# B&R Automation Studio project testovaci_pneu_stan (part 2)

#### regulatory.fun
```iecst
FUNCTION_BLOCK FF_PID_r_t
	VAR_INPUT
		ssMethodType :  SINT;
		stiffness_ff :  REAL :=  0; (*tuhos ff regulatora (sum tlakov)*)
		ref_alfa_x :  REAL :=  0; (*requested alfa x in deg*)
		ref_alfa_y :  REAL :=  0; (*requested alfa y in deg*)
		real_alfa_x :  REAL :=  0; (*requested alfa x in deg*)
		real_alfa_y :  REAL :=  0; (*requested alfa y in deg*)
		P_parameter :  REAL :=  0; (*parameter P PID*)
		reset_PID_blue :  REAL :=  0; (*requested alfa x in deg*)
		D_parameter :  REAL :=  0; (*parameter D PID*)
		N_parameter :  REAL :=  0; (*parameter N PID*)
		reset_PID_green :  REAL :=  0; (*requested alfa x in deg*)
		reset_PID_yellow :  REAL :=  0; (*requested alfa x in deg*)
		tlak3 :  REAL :=  0; (*aktu&#xFFFD; (*aktu&#xFFFD;lny tlak green*)
		I_parameter :  REAL :=  0; (*parameter I PID*)
		tlak1 :  REAL :=  0; (*aktu&#xFFFD; (*aktu&#xFFFD;lny tlak blue*)
		tlak2 :  REAL :=  0; (*aktu&#xFFFD; (*aktu&#xFFFD;lny tlak yellow*)
	END_VAR
	VAR_OUTPUT
		Blue_tab :  REAL :=  0; (*Blue_pressure*)
		Yellow_tab :  REAL :=  0; (*Yellow_pressure*)
		Green_tab :  REAL :=  0; (*Green_pressure*)
	END_VAR
	VAR
		bur_B_reg_FF_PI_pl_regr_stiff_T :  B_reg_FF_PI_pl_regr_stiff_T;
		bur_DW_reg_FF_PI_pl_regr_stiff_ :  DW_reg_FF_PI_pl_regr_stiff_T;
		bur_reg_FF_PI_pl_regr_stiff :  tag_RTM_reg_FF_PI_pl_regr_sti_T;
	END_VAR
END_FUNCTION_BLOCK

FUNCTION_BLOCK PID_c
	VAR_INPUT
		ssMethodType :  SINT;
		ref_alfa_x :  REAL :=   0; (*requested alfa x in deg*)
		ref_alfa_y :  REAL :=   0; (*requested alfa y in deg*)
		real_alfa_x :  REAL :=   0; (*requested alfa x in deg*)
		real_alfa_y :  REAL :=   0; (*requested alfa y in deg*)
		P_parameter :  REAL :=   0; (*parameter P PID*)
		reset_PID_blue :  REAL :=   0; (*requested alfa x in deg*)
		D_parameter :  REAL :=   0; (*parameter D PID*)
		N_parameter :  REAL :=   0; (*parameter N PID*)
		reset_PID_yellow :  REAL :=   0; (*requested alfa x in deg*)
		reset_PID_green :  REAL :=   0; (*requested alfa x in deg*)
		I_parameter :  REAL :=   0; (*parameter I PID*)
	END_VAR
	VAR_OUTPUT
		Blue_tab :  REAL :=   0; (*Blue_pressure*)
		Yellow_tab :  REAL :=   0; (*Yellow_pressure*)
		Green_tab :  REAL :=   0; (*Green_pressure*)
	END_VAR
	VAR
		bur_B_PID_co_T :  B_PID_co_T;
		bur_DW_PID_co_T :  DW_PID_co_T;
		bur_PID_co :  tag_RTM_PID_co_T;
	END_VAR
END_FUNCTION_BLOCK

FUNCTION_BLOCK nonL_P
	VAR_INPUT
		ssMethodType :  SINT;
		ref_alfa_x :  REAL :=     0; (*requested alfa x in deg*)
		ref_alfa_y :  REAL :=     0; (*requested alfa y in deg*)
		real_alfa_x :  REAL :=     0; (*requested alfa x in deg*)
		real_alfa_y :  REAL :=     0; (*requested alfa y in deg*)
	END_VAR
	VAR_OUTPUT
		Blue_tab :  REAL :=     0; (*Blue_pressure*)
		Yellow_tab :  REAL :=     0; (*Yellow_pressure*)
		Green_tab :  REAL :=     0; (*Green_pressure*)
	END_VAR
	VAR
		bur_B_regulator_nelin_P_T :  B_regulator_nelin_P_T;
		bur_regulator_nelin_P :  tag_RTM_regulator_nelin_P_T;
	END_VAR
END_FUNCTION_BLOCK

FUNCTION_BLOCK FF_PID_r
	VAR_INPUT
		ssMethodType :  SINT;
		ref_alfa_x :  REAL :=         0; (*requested alfa x in deg*)
		ref_alfa_y :  REAL :=         0; (*requested alfa y in deg*)
		real_alfa_x :  REAL :=         0; (*requested alfa x in deg*)
		real_alfa_y :  REAL :=         0; (*requested alfa y in deg*)
		P_parameter :  REAL :=         0; (*parameter P PID*)
		reset_PID_blue :  REAL :=         0; (*requested alfa x in deg*)
		D_parameter :  REAL :=         0; (*parameter D PID*)
		N_parameter :  REAL :=         0; (*parameter N PID*)
		reset_PID_green :  REAL :=         0; (*requested alfa x in deg*)
		reset_PID_yellow :  REAL :=         0; (*requested alfa x in deg*)
		tlak3 :  REAL :=         0; (*aktu&#xFFFD; (*aktu&#xFFFD; (*aktu&#xFFFD; (*aktu&#xFFFD; (*aktu&#xFFFD; (*aktu&#xFFFD; (*aktu&#xFFFD; (*aktu&#xFFFD; (*aktu&#xFFFD; (*aktu&#xFFFD; (*aktu&#xFFFD; (*aktu&#xFFFD; (*aktu&#xFFFD; (*aktu&#xFFFD; (*aktu&#xFFFD; (*aktu&#xFFFD; (*aktu&#xFFFD; (*aktu&#xFFFD; (*aktu&#xFFFD; (*aktu&#xFFFD; (*aktu&#xFFFD; (*aktu&#xFFFD; (*aktu&#xFFFD; (*aktu&#xFFFD; (*aktu&#xFFFD; (*aktu&#xFFFD; (*aktu&#xFFFD; (*aktu&#xFFFD; (*aktu&#xFFFD; (*aktu&#xFFFD; (*aktu&#xFFFD; (*aktu&#xFFFD; (*aktu&#xFFFD; (*aktu&#xFFFD; (*aktu&#xFFFD; (*aktu&#xFFFD; (*aktu&#xFFFD; (*aktu&#xFFFD; (*aktu&#xFFFD; (*aktu&#xFFFD; (*aktu&#xFFFD; (*aktu&#xFFFD; (*aktu&#xFFFD; (*aktu&#xFFFD; (*aktu&#xFFFD; (*aktu&#xFFFD; (*aktu&#xFFFD; (*aktu&#xFFFD; (*aktu&#xFFFD; (*aktu&#xFFFD; (*aktu&#xFFFD; (*aktu&#xFFFD; (*aktu&#xFFFD; (*aktu&#xFFFD; (*aktu&#xFFFD; (*aktu&#xFFFD; (*aktu&#xFFFD; (*aktu&#xFFFD; (*aktu&#xFFFD; (*aktu&#xFFFD; (*aktu&#xFFFD; (*aktu&#xFFFD; (*aktu&#xFFFD; (*aktu&#xFFFD; (*aktu&#xFFFD; (*aktu&#xFFFD; (*aktu&#xFFFD; (*aktu&#xFFFD; (*aktu&#xFFFD; (*aktu&#xFFFD; (*aktu&#xFFFD; (*aktu&#xFFFD; (*aktu&#xFFFD; (*aktu&#xFFFD; (*aktu&#xFFFD; (*aktu&#xFFFD; (*aktu&#xFFFD; (*aktu&#xFFFD; (*aktu&#xFFFD; (*aktu&#xFFFD; (*aktu&#xFFFD; (*aktu&#xFFFD; (*aktu&#xFFFD; (*aktu&#xFFFD; (*aktu&#xFFFD; (*aktu&#xFFFD; (*aktu&#xFFFD; (*aktu&#xFFFD; (*aktu&#xFFFD; (*aktu&#xFFFD; (*aktu&#xFFFD; (*aktu&#xFFFD; (*aktu&#xFFFD; (*aktu&#xFFFD; (*aktu&#xFFFD; (*aktu&#xFFFD; (*aktu&#xFFFD; (*aktu&#xFFFD; (*aktu&#xFFFD; (*aktu&#xFFFD; (*aktu&#xFFFD; (*aktu&#xFFFD; (*aktu&#xFFFD; (*aktu&#xFFFD; (*aktu&#xFFFD; (*aktu&#xFFFD; (*aktu&#xFFFD; (*aktu&#xFFFD; (*aktu&#xFFFD; (*aktu&#xFFFD; (*aktu&#xFFFD; (*aktu&#xFFFD; (*aktu&#xFFFD; (*aktu&#xFFFD; (*aktu&#xFFFD; (*aktu&#xFFFD; (*aktu&#xFFFD; (*aktu&#xFFFD; (*aktu&#xFFFD; (*aktu&#xFFFD; (*aktu&#xFFFD; (*aktu&#xFFFD; (*aktu&#xFFFD; (*aktu&#xFFFD; (*aktu&#xFFFD; (*aktu&#xFFFD; (*aktu&#xFFFD; (*aktu&#xFFFD; (*aktu&#xFFFD; (*aktu&#xFFFD; (*aktu&#xFFFD; (*aktu&#xFFFD; (*aktu&#xFFFD; (*aktu&#xFFFD; (*aktu&#xFFFD; (*aktu&#xFFFD; (*aktu&#xFFFD; (*aktu&#xFFFD; (*aktu&#xFFFD; (*aktu&#xFFFD; (*aktu&#xFFFD; (*aktu&#xFFFD; (*aktu&#xFFFD; (*aktu&#xFFFD; (*aktu&#xFFFD; (*aktu&#xFFFD; (*aktu&#xFFFD; (*aktu&#xFFFD; (*aktu&#xFFFD; (*aktu&#xFFFD; (*aktu&#xFFFD; (*aktu&#xFFFD; (*aktu&#xFFFD; (*aktu&#xFFFD; (*aktu&#xFFFD; (*aktu&#xFFFD; (*aktu&#xFFFD; (*aktu&#xFFFD; (*aktu&#xFFFD; (*aktu&#xFFFD; (*aktu&#xFFFD; (*aktu&#xFFFD; (*aktu&#xFFFD; (*aktu&#xFFFD; (*aktu&#xFFFD; (*aktu&#xFFFD; (*aktu&#xFFFD; (*aktu&#xFFFD; (*aktu&#xFFFD; (*aktu&#xFFFD; (*aktu&#xFFFD; (*aktu&#xFFFD; (*aktu&#xFFFD; (*aktu&#xFFFD; (*aktu&#xFFFD; (*aktu&#xFFFD; (*aktu&#xFFFD; (*aktu&#xFFFD; (*aktu&#xFFFD; (*aktu&#xFFFD; (*aktu&#xFFFD; (*aktu&#xFFFD; (*aktu&#xFFFD; (*aktu&#xFFFD; (*aktu&#xFFFD; (*aktu&#xFFFD; (*aktu&#xFFFD; (*aktu&#xFFFD; (*aktu&#xFFFD; (*aktu&#xFFFD; (*aktu&#xFFFD; (*aktu&#xFFFD; (*aktu&#xFFFD; (*aktu&#xFFFD; (*aktu&#xFFFD; (*aktu&#xFFFD; (*aktu&#xFFFD; (*aktu&#xFFFD; (*aktu&#xFFFD; (*aktu&#xFFFD; (*aktu&#xFFFD; (*aktu&#xFFFD; (*aktu&#xFFFD; (*aktu&#xFFFD; (*aktu&#xFFFD; (*aktu&#xFFFD; (*aktu&#xFFFD; (*aktu&#xFFFD; (*aktu&#xFFFD; (*aktu&#xFFFD; (*aktu&#xFFFD; (*aktu&#xFFFD; (*aktu&#xFFFD; (*aktu&#xFFFD; (*aktu&#xFFFD; (*aktu&#xFFFD; (*aktu&#xFFFD; (*aktu&#xFFFD; (*aktu&#xFFFD; (*aktu&#xFFFD; (*aktu&#xFFFD; (*aktu&#xFFFD; (*aktu&#xFFFD; (*aktu&#xFFFD; (*aktu&#xFFFD; (*aktu&#xFFFD; (*aktu&#xFFFD; (*aktu&#xFFFD; (*aktu&#xFFFD; (*aktu&#xFFFD; (*aktu&#xFFFD; (*aktu&#xFFFD; (*aktu&#xFFFD; (*aktu&#xFFFD; (*aktu&#xFFFD; (*aktu&#xFFFD; (*aktu&#xFFFD; (*aktu&#xFFFD; (*aktu&#xFFFD; (*aktu&#xFFFD; (*aktu&#xFFFD; (*aktu&#xFFFD; (*aktu&#xFFFD; (*aktu&#xFFFD; (*aktu&#xFFFD; (*aktu&#xFFFD; (*aktu&#xFFFD; (*aktu&#xFFFD; (*aktu&#xFFFD; (*aktu&#xFFFD; (*aktu&#xFFFD; (*aktu&#xFFFD; (*aktu&#xFFFD; (*aktu&#xFFFD; (*aktu&#xFFFD; (*aktu&#xFFFD; (*aktu&#xFFFD; (*aktu&#xFFFD; (*aktu&#xFFFD; (*aktu&#xFFFD; (*aktu&#xFFFD; (*aktu&#xFFFD; (*aktu&#xFFFD; (*aktu&#xFFFD; (*aktu&#xFFFD; (*aktu&#xFFFD; (*aktu&#xFFFD; (*aktu&#xFFFD; (*aktu&#xFFFD; (*aktu&#xFFFD; (*aktu&#xFFFD; (*aktu&#xFFFD; (*aktu&#xFFFD; (*aktu&#xFFFD; (*aktu&#xFFFD; (*aktu&#xFFFD; (*aktu&#xFFFD; (*aktu&#xFFFD; (*aktu&#xFFFD; (*aktu&#xFFFD; (*aktu&#xFFFD; (*aktu&#xFFFD; (*aktu&#xFFFD; (*aktu&#xFFFD; (*aktu&#xFFFD; (*aktu&#xFFFD; (*aktu&#xFFFD; (*aktu&#xFFFD; (*aktu&#xFFFD; (*aktu&#xFFFD; (*aktu&#xFFFD; (*aktu&#xFFFD; (*aktu&#xFFFD; (*aktu&#xFFFD; (*aktu&#xFFFD; (*aktu&#xFFFD; (*aktu&#xFFFD; (*aktu&#xFFFD; (*aktu&#xFFFD; (*aktu&#xFFFD; (*aktu&#xFFFD; (*aktu&#xFFFD; (*aktu&#xFFFD; (*aktu&#xFFFD; (*aktu&#xFFFD; (*aktu&#xFFFD; (*aktu&#xFFFD; (*aktu&#xFFFD; (*aktu&#xFFFD; (*aktu&#xFFFD; (*aktu&#xFFFD; (*aktu&#xFFFD; (*aktu&#xFFFD; (*aktu&#xFFFD; (*aktu&#xFFFD; (*aktu&#xFFFD; (*aktu&#xFFFD; (*aktu&#xFFFD; (*aktu&#xFFFD; (*aktu&#xFFFD; (*aktu&#xFFFD; (*aktu&#xFFFD; (*aktu&#xFFFD; (*aktu&#xFFFD; (*aktu&#xFFFD; (*aktu&#xFFFD; (*aktu&#xFFFD; (*aktu&#xFFFD; (*aktu&#xFFFD; (*aktu&#xFFFD; (*aktu&#xFFFD; (*aktu&#xFFFD; (*aktu&#xFFFD; (*aktu&#xFFFD; (*aktu&#xFFFD; (*aktu&#xFFFD; (*aktu&#xFFFD; (*aktu&#xFFFD; (*aktu&#xFFFD; (*aktu&#xFFFD; (*aktu&#xFFFD; (*aktu&#xFFFD; (*aktu&#xFFFD; (*aktu&#xFFFD; (*aktu&#xFFFD; (*aktu&#xFFFD; (*aktu&#xFFFD; (*aktu&#xFFFD; (*aktu&#xFFFD; (*aktu&#xFFFD; (*aktu&#xFFFD; (*aktu&#xFFFD; (*aktu&#xFFFD; (*aktu&#xFFFD; (*aktu&#xFFFD; (*aktu&#xFFFD; (*aktu&#xFFFD; (*aktu&#xFFFD; (*aktu&#xFFFD; (*aktu&#xFFFD; (*aktu&#xFFFD; (*aktu&#xFFFD; (*aktu&#xFFFD; (*aktu&#xFFFD; (*aktu&#xFFFD; (*aktu&#xFFFD; (*aktu&#xFFFD; (*aktu&#xFFFD; (*aktu&#xFFFD; (*aktu&#xFFFD; (*aktu&#xFFFD; (*aktu&#xFFFD; (*aktu&#xFFFD; (*aktu&#xFFFD; (*aktu&#xFFFD; (*aktu&#xFFFD; (*aktu&#xFFFD; (*aktu&#xFFFD; (*aktu&#xFFFD; (*aktu&#xFFFD; (*aktu&#xFFFD; (*aktu&#xFFFD; (*aktu&#xFFFD; (*aktu&#xFFFD; (*aktu&#xFFFD; (*aktu&#xFFFD; (*aktu&#xFFFD; (*aktu&#xFFFD; (*aktu&#xFFFD; (*aktu&#xFFFD; (*aktu&#xFFFD; (*aktu&#xFFFD; (*aktu&#xFFFD; (*aktu&#xFFFD; (*aktu&#xFFFD; (*aktu&#xFFFD; (*aktu&#xFFFD; (*aktu&#xFFFD; (*aktu&#xFFFD; (*aktu&#xFFFD; (*aktu&#xFFFD; (*aktu&#xFFFD; (*aktu&#xFFFD; (*aktu&#xFFFD; (*aktu&#xFFFD; (*aktu&#xFFFD; (*aktu&#xFFFD; (*aktu&#xFFFD; (*aktu&#xFFFD; (*aktu&#xFFFD; (*aktu&#xFFFD; (*aktu&#xFFFD; (*aktu&#xFFFD; (*aktu&#xFFFD; (*aktu&#xFFFD; (*aktu&#xFFFD; (*aktu&#xFFFD; (*aktu&#xFFFD; (*aktu&#xFFFD; (*aktu&#xFFFD; (*aktu&#xFFFD; (*aktu&#xFFFD; (*aktu&#xFFFD; (*aktu&#xFFFD; (*aktu&#xFFFD; (*aktu&#xFFFD; (*aktu&#xFFFD; (*aktu&#xFFFD; (*aktu&#xFFFD; (*aktu&#xFFFD; (*aktu&#xFFFD; (*aktu&#xFFFD; (*aktu&#xFFFD; (*aktu&#xFFFD; (*aktu&#xFFFD; (*aktu&#xFFFD; (*aktu&#xFFFD; (*aktu&#xFFFD; (*aktu&#xFFFD; (*aktu&#xFFFD; (*aktu&#xFFFD; (*aktu&#xFFFD; (*aktu&#xFFFD; (*aktu&#xFFFD; (*aktu&#xFFFD; (*aktu&#xFFFD; (*aktu&#xFFFD; (*aktu&#xFFFD; (*aktu&#xFFFD; (*aktu&#xFFFD; (*aktu&#xFFFD; (*aktu&#xFFFD; (*aktu&#xFFFD; (*aktu&#xFFFD; (*aktu&#xFFFD; (*aktu&#xFFFD; (*aktu&#xFFFD; (*aktu&#xFFFD; (*aktu&#xFFFD; (*aktu&#xFFFD; (*aktu&#xFFFD; (*aktu&#xFFFD; (*aktu&#xFFFD; (*aktu&#xFFFD; (*aktu&#xFFFD; (*aktu&#xFFFD; (*aktu&#xFFFD; (*aktu&#xFFFD; (*aktu&#xFFFD; (*aktu&#xFFFD; (*aktu&#xFFFD; (*aktu&#xFFFD; (*aktu&#xFFFD; (*aktu&#xFFFD; (*aktu&#xFFFD; (*aktu&#xFFFD; (*aktu&#xFFFD; (*aktu&#xFFFD; (*aktu&#xFFFD; (*aktu&#xFFFD; (*aktu&#xFFFD; (*aktu&#xFFFD; (*aktu&#xFFFD; (*aktu&#xFFFD; (*aktu&#xFFFD; (*aktu&#xFFFD; (*aktu&#xFFFD; (*aktu&#xFFFD; (*aktu&#xFFFD; (*aktu&#xFFFD; (*aktu&#xFFFD; (*aktu&#xFFFD; (*aktu&#xFFFD; (*aktu&#xFFFD; (*aktu&#xFFFD; (*aktu&#xFFFD; (*aktu&#xFFFD; (*aktu&#xFFFD; (*aktu&#xFFFD; (*aktu&#xFFFD; (*aktu&#xFFFD; (*aktu&#xFFFD; (*aktu&#xFFFD; (*aktu&#xFFFD; (*aktu&#xFFFD; (*aktu&#xFFFD; (*aktu&#xFFFD; (*aktu&#xFFFD; (*aktu&#xFFFD; (*aktu&#xFFFD; (*aktu&#xFFFD; (*aktu&#xFFFD; (*aktu&#xFFFD; (*aktu&#xFFFD; (*aktu&#xFFFD; (*aktu&#xFFFD; (*aktu&#xFFFD; (*aktu&#xFFFD; (*aktu&#xFFFD; (*aktu&#xFFFD; (*aktu&#xFFFD; (*aktu&#xFFFD; (*aktu&#xFFFD; (*aktu&#xFFFD; (*aktu&#xFFFD; (*aktu&#xFFFD; (*aktu&#xFFFD; (*aktu&#xFFFD; (*aktu&#xFFFD; (*aktu&#xFFFD; (*aktu&#xFFFD; (*aktu&#xFFFD; (*aktu&#xFFFD; (*aktu&#xFFFD; (*aktu&#xFFFD; (*aktu&#xFFFD; (*aktu&#xFFFD; (*aktu&#xFFFD; (*aktu&#xFFFD; (*aktu&#xFFFD; (*aktu&#xFFFD; (*aktu&#xFFFD; (*aktu&#xFFFD; (*aktu&#xFFFD; (*aktu&#xFFFD; (*aktu&#xFFFD; (*aktu&#xFFFD; (*aktu&#xFFFD; (*aktu&#xFFFD; (*aktu&#xFFFD; (*aktu&#xFFFD; (*aktu&#xFFFD; (*aktu&#xFFFD; (*aktu&#xFFFD; (*aktu&#xFFFD; (*aktu&#xFFFD; (*aktu&#xFFFD; (*aktu&#xFFFD; (*aktu&#xFFFD; (*aktu&#xFFFD; (*aktu&#xFFFD; (*aktu&#xFFFD; (*aktu&#xFFFD; (*aktu&#xFFFD; (*aktu&#xFFFD; (*aktu&#xFFFD; (*aktu&#xFFFD; (*aktu&#xFFFD; (*aktu&#xFFFD; (*aktu&#xFFFD; (*aktu&#xFFFD; (*aktu&#xFFFD; (*aktu&#xFFFD; (*aktu&#xFFFD; (*aktu&#xFFFD; (*aktu&#xFFFD; (*aktu&#xFFFD; (*aktu&#xFFFD; (*aktu&#xFFFD; (*aktu&#xFFFD; (*aktu&#xFFFD; (*aktu&#xFFFD; (*aktu&#xFFFD; (*aktu&#xFFFD; (*aktu&#xFFFD; (*aktu&#xFFFD; (*aktu&#xFFFD; (*aktu&#xFFFD; (*aktu&#xFFFD; (*aktu&#xFFFD; (*aktu&#xFFFD; (*aktu&#xFFFD; (*aktu&#xFFFD; (*aktu&#xFFFD; (*aktu&#xFFFD; (*aktu&#xFFFD; (*aktu&#xFFFD; (*aktu&#xFFFD; (*aktu&#xFFFD; (*aktu&#xFFFD; (*aktu&#xFFFD; (*aktu&#xFFFD; (*aktu&#xFFFD; (*aktu&#xFFFD; (*aktu&#xFFFD; (*aktu&#xFFFD; (*aktu&#xFFFD; (*aktu&#xFFFD; (*aktu&#xFFFD; (*aktu&#xFFFD; (*aktu&#xFFFD; (*aktu&#xFFFD; (*aktu&#xFFFD; (*aktu&#xFFFD; (*aktu&#xFFFD; (*aktu&#xFFFD; (*aktu&#xFFFD; (*aktu&#xFFFD; (*aktu&#xFFFD; (*aktu&#xFFFD; (*aktu&#xFFFD; (*aktu&#xFFFD; (*aktu&#xFFFD; (*aktu&#xFFFD; (*aktu&#xFFFD; (*aktu&#xFFFD; (*aktu&#xFFFD; (*aktu&#xFFFD; (*aktu&#xFFFD; (*aktu&#xFFFD; (*aktu&#xFFFD; (*aktu&#xFFFD; (*aktu&#xFFFD; (*aktu&#xFFFD; (*aktu&#xFFFD; (*aktu&#xFFFD; (*aktu&#xFFFD; (*aktu&#xFFFD; (*aktu&#xFFFD; (*aktu&#xFFFD; (*aktu&#xFFFD; (*aktu&#xFFFD; (*aktu&#xFFFD; (*aktu&#xFFFD; (*aktu&#xFFFD; (*aktu&#xFFFD; (*aktu&#xFFFD; (*aktu&#xFFFD; (*aktu&#xFFFD; (*aktu&#xFFFD; (*aktu&#xFFFD; (*aktu&#xFFFD; (*aktu&#xFFFD; (*aktu&#xFFFD; (*aktu&#xFFFD; (*aktu&#xFFFD; (*aktu&#xFFFD; (*aktu&#xFFFD; (*aktu&#xFFFD; (*aktu&#xFFFD; (*aktu&#xFFFD; (*aktu&#xFFFD; (*aktu&#xFFFD; (*aktu&#xFFFD; (*aktu&#xFFFD; (*aktu&#xFFFD; (*aktu&#xFFFD; (*aktu&#xFFFD; (*aktu&#xFFFD; (*aktu&#xFFFD; (*aktu&#xFFFD; (*aktu&#xFFFD; (*aktu&#xFFFD; (*aktu&#xFFFD; (*aktu&#xFFFD; (*aktu&#xFFFD; (*aktu&#xFFFD; (*aktu&#xFFFD; (*aktu&#xFFFD; (*aktu&#xFFFD; (*aktu&#xFFFD; (*aktu&#xFFFD; (*aktu&#xFFFD; (*aktu&#xFFFD; (*aktu&#xFFFD; (*aktu&#xFFFD; (*aktu&#xFFFD; (*aktu&#xFFFD; (*aktu&#xFFFD; (*aktu&#xFFFD; (*aktu&#xFFFD; (*aktu&#xFFFD; (*aktu&#xFFFD; (*aktu&#xFFFD; (*aktu&#xFFFD; (*aktu&#xFFFD; (*aktu&#xFFFD; (*aktu&#xFFFD; (*aktu&#xFFFD; (*aktu&#xFFFD; (*aktu&#xFFFD; (*aktu&#xFFFD; (*aktu&#xFFFD; (*aktu&#xFFFD; (*aktu&#xFFFD; (*aktu&#xFFFD; (*aktu&#xFFFD; (*aktu&#xFFFD; (*aktu&#xFFFD; (*aktu&#xFFFD; (*aktu&#xFFFD; (*aktu&#xFFFD; (*aktu&#xFFFD; (*aktu&#xFFFD; (*aktu&#xFFFD; (*aktu&#xFFFD; (*aktu&#xFFFD; (*aktu&#xFFFD; (*aktu&#xFFFD; (*aktu&#xFFFD; (*aktu&#xFFFD; (*aktu&#xFFFD; (*aktu&#xFFFD; (*aktu&#xFFFD; (*aktu&#xFFFD; (*aktu&#xFFFD; (*aktu&#xFFFD; (*aktu&#xFFFD; (*aktu&#xFFFD; (*aktu&#xFFFD; (*aktu&#xFFFD; (*aktu&#xFFFD; (*aktu&#xFFFD; (*aktu&#xFFFD; (*aktu&#xFFFD; (*aktu&#xFFFD; (*aktu&#xFFFD; (*aktu&#xFFFD; (*aktu&#xFFFD; (*aktu&#xFFFD; (*aktu&#xFFFD; (*aktu&#xFFFD; (*aktu&#xFFFD; (*aktu&#xFFFD; (*aktu&#xFFFD; (*aktu&#xFFFD; (*aktu&#xFFFD; (*aktu&#xFFFD; (*aktu&#xFFFD; (*aktu&#xFFFD; (*aktu&#xFFFD; (*aktu&#xFFFD; (*aktu&#xFFFD; (*aktu&#xFFFD; (*aktu&#xFFFD; (*aktu&#xFFFD; (*aktu&#xFFFD; (*aktu&#xFFFD; (*aktu&#xFFFD; (*aktu&#xFFFD; (*aktu&#xFFFD; (*aktu&#xFFFD; (*aktu&#xFFFD; (*aktu&#xFFFD; (*aktu&#xFFFD; (*aktu&#xFFFD; (*aktu&#xFFFD; (*aktu&#xFFFD; (*aktu&#xFFFD; (*aktu&#xFFFD; (*aktu&#xFFFD; (*aktu&#xFFFD; (*aktu&#xFFFD; (*aktu&#xFFFD; (*aktu&#xFFFD; (*aktu&#xFFFD; (*aktu&#xFFFD; (*aktu&#xFFFD; (*aktu&#xFFFD; (*aktu&#xFFFD; (*aktu&#xFFFD; (*aktu&#xFFFD; (*aktu&#xFFFD; (*aktu&#xFFFD; (*aktu&#xFFFD; (*aktu&#xFFFD; (*aktu&#xFFFD; (*aktu&#xFFFD; (*aktu&#xFFFD; (*aktu&#xFFFD; (*aktu&#xFFFD; (*aktu&#xFFFD; (*aktu&#xFFFD; (*aktu&#xFFFD; (*aktu&#xFFFD; (*aktu&#xFFFD; (*aktu&#xFFFD; (*aktu&#xFFFD; (*aktu&#xFFFD; (*aktu&#xFFFD; (*aktu&#xFFFD; (*aktu&#xFFFD; (*aktu&#xFFFD; (*aktu&#xFFFD; (*aktu&#xFFFD; (*aktu&#xFFFD; (*aktu&#xFFFD; (*aktu&#xFFFD; (*aktu&#xFFFD; (*aktu&#xFFFD; (*aktu&#xFFFD; (*aktu&#xFFFD; (*aktu&#xFFFD; (*aktu&#xFFFD; (*aktu&#xFFFD; (*aktu&#xFFFD; (*aktu&#xFFFD; (*aktu&#xFFFD; (*aktu&#xFFFD; (*aktu&#xFFFD; (*aktu&#xFFFD; (*aktu&#xFFFD; (*aktu&#xFFFD; (*aktu&#xFFFD; (*aktu&#xFFFD; (*aktu&#xFFFD; (*aktu&#xFFFD; (*aktu&#xFFFD; (*aktu&#xFFFD; (*aktu&#xFFFD; (*aktu&#xFFFD; (*aktu&#xFFFD; (*aktu&#xFFFD; (*aktu&#xFFFD; (*aktu&#xFFFD; (*aktu&#xFFFD; (*aktu&#xFFFD; (*aktu&#xFFFD; (*aktu&#xFFFD; (*aktu&#xFFFD; (*aktu&#xFFFD; (*aktu&#xFFFD; (*aktu&#xFFFD; (*aktu&#xFFFD; (*aktu&#xFFFD; (*aktu&#xFFFD; (*aktu&#xFFFD; (*aktu&#xFFFD; (*aktu&#xFFFD; (*aktu&#xFFFD; (*aktu&#xFFFD; (*aktu&#xFFFD; (*aktu&#xFFFD; (*aktu&#xFFFD; (*aktu&#xFFFD; (*aktu&#xFFFD; (*aktu&#xFFFD; (*aktu&#xFFFD; (*aktu&#xFFFD; (*aktu&#xFFFD; (*aktu&#xFFFD; (*aktu&#xFFFD; (*aktu&#xFFFD; (*aktu&#xFFFD; (*aktu&#xFFFD; (*aktu&#xFFFD; (*aktu&#xFFFD; (*aktu&#xFFFD; (*aktu&#xFFFD; (*aktu&#xFFFD; (*aktu&#xFFFD; (*aktu&#xFFFD; (*aktu&#xFFFD; (*aktu&#xFFFD; (*aktu&#xFFFD; (*aktu&#xFFFD; (*aktu&#xFFFD; (*aktu&#xFFFD; (*aktu&#xFFFD; (*aktu&#xFFFD; (*aktu&#xFFFD; (*aktu&#xFFFD; (*aktu&#xFFFD; (*aktu&#xFFFD; (*aktu&#xFFFD; (*aktu&#xFFFD; (*aktu&#xFFFD; (*aktu&#xFFFD; (*aktu&#xFFFD; (*aktu&#xFFFD; (*aktu&#xFFFD; (*aktu&#xFFFD; (*aktu&#xFFFD; (*aktu&#xFFFD; (*aktu&#xFFFD; (*aktu&#xFFFD; (*aktu&#xFFFD; (*aktu&#xFFFD; (*aktu&#xFFFD; (*aktu&#xFFFD; (*aktu&#xFFFD; (*aktu&#xFFFD; (*aktu&#xFFFD; (*aktu&#xFFFD; (*aktu&#xFFFD; (*aktu&#xFFFD; (*aktu&#xFFFD; (*aktu&#xFFFD; (*aktu&#xFFFD; (*aktu&#xFFFD; (*aktu&#xFFFD; (*aktu&#xFFFD; (*aktu&#xFFFD; (*aktu&#xFFFD; (*aktu&#xFFFD; (*aktu&#xFFFD; (*aktu&#xFFFD; (*aktu&#xFFFD; (*aktu&#xFFFD; (*aktu&#xFFFD; (*aktu&#xFFFD; (*aktu&#xFFFD; (*aktu&#xFFFD; (*aktu&#xFFFD; (*aktu&#xFFFD; (*aktu&#xFFFD; (*aktu&#xFFFD; (*aktu&#xFFFD; (*aktu&#xFFFD; (*aktu&#xFFFD; (*aktu&#xFFFD; (*aktu&#xFFFD; (*aktu&#xFFFD; (*aktu&#xFFFD; (*aktu&#xFFFD; (*aktu&#xFFFD; (*aktu&#xFFFD; (*aktu&#xFFFD; (*aktu&#xFFFD; (*aktu&#xFFFD; (*aktu&#xFFFD; (*aktu&#xFFFD; (*aktu&#xFFFD; (*aktu&#xFFFD; (*aktu&#xFFFD; (*aktu&#xFFFD; (*aktu&#xFFFD; (*aktu&#xFFFD; (*aktu&#xFFFD; (*aktu&#xFFFD; (*aktu&#xFFFD; (*aktu&#xFFFD; (*aktu&#xFFFD; (*aktu&#xFFFD; (*aktu&#xFFFD; (*aktu&#xFFFD; (*aktu&#xFFFD; (*aktu&#xFFFD; (*aktu&#xFFFD; (*aktu&#xFFFD; (*aktu&#xFFFD; (*aktu&#xFFFD; (*aktu&#xFFFD; (*aktu&#xFFFD; (*aktu&#xFFFD; (*aktu&#xFFFD; (*aktu&#xFFFD; (*aktu&#xFFFD; (*aktu&#xFFFD; (*aktu&#xFFFD; (*aktu&#xFFFD; (*aktu&#xFFFD; (*aktu&#xFFFD; (*aktu&#xFFFD; (*aktu&#xFFFD; (*aktu&#xFFFD; (*aktu&#xFFFD; (*aktu&#xFFFD; (*aktu&#xFFFD; (*aktu&#xFFFD; (*aktu&#xFFFD; (*aktu&#xFFFD; (*aktu&#xFFFD; (*aktu&#xFFFD; (*aktu&#xFFFD; (*aktu&#xFFFD; (*aktu&#xFFFD; (*aktu&#xFFFD; (*aktu&#xFFFD; (*aktu&#xFFFD; (*aktu&#xFFFD; (*aktu&#xFFFD; (*aktu&#xFFFD; (*aktu&#xFFFD; (*aktu&#xFFFD; (*aktu&#xFFFD; (*aktu&#xFFFD; (*aktu&#xFFFD; (*aktu&#xFFFD; (*aktu&#xFFFD; (*aktu&#xFFFD; (*aktu&#xFFFD; (*aktu&#xFFFD; (*aktu&#xFFFD; (*aktu&#xFFFD; (*aktu&#xFFFD; (*aktu&#xFFFD; (*aktu&#xFFFD; (*aktu&#xFFFD; (*aktu&#xFFFD; (*aktu&#xFFFD; (*aktu&#xFFFD; (*aktu&#xFFFD; (*aktu&#xFFFD; (*aktu&#xFFFD; (*aktu&#xFFFD; (*aktu&#xFFFD; (*aktu&#xFFFD; (*aktu&#xFFFD; (*aktu&#xFFFD; (*aktu&#xFFFD; (*aktu&#xFFFD; (*aktu&#xFFFD; (*aktu&#xFFFD; (*aktu&#xFFFD; (*aktu&#xFFFD; (*aktu&#xFFFD; (*aktu&#xFFFD; (*aktu&#xFFFD; (*aktu&#xFFFD; (*aktu&#xFFFD; (*aktu&#xFFFD; (*aktu&#xFFFD; (*aktu&#xFFFD; (*aktu&#xFFFD; (*aktu&#xFFFD; (*aktu&#xFFFD; (*aktu&#xFFFD; (*aktu&#xFFFD; (*aktu&#xFFFD; (*aktu&#xFFFD; (*aktu&#xFFFD; (*aktu&#xFFFD; (*aktu&#xFFFD; (*aktu&#xFFFD; (*aktu&#xFFFD; (*aktu&#xFFFD; (*aktu&#xFFFD; (*aktu&#xFFFD; (*aktu&#xFFFD; (*aktu&#xFFFD; (*aktu&#xFFFD; (*aktu&#xFFFD; (*aktu&#xFFFD; (*aktu&#xFFFD; (*aktu&#xFFFD; (*aktu&#xFFFD; (*aktu&#xFFFD; (*aktu&#xFFFD; (*aktu&#xFFFD; (*aktu&#xFFFD; (*aktu&#xFFFD; (*aktu&#xFFFD; (*aktu&#xFFFD; (*aktu&#xFFFD; (*aktu&#xFFFD; (*aktu&#xFFFD; (*aktu&#xFFFD; (*aktu&#xFFFD; (*aktu&#xFFFD; (*aktu&#xFFFD; (*aktu&#xFFFD; (*aktu&#xFFFD; (*aktu&#xFFFD; (*aktu&#xFFFD; (*aktu&#xFFFD; (*aktu&#xFFFD; (*aktu&#xFFFD; (*aktu&#xFFFD; (*aktu&#xFFFD; (*aktu&#xFFFD; (*aktu&#xFFFD; (*aktu&#xFFFD; (*aktu&#xFFFD; (*aktu&#xFFFD; (*aktu&#xFFFD; (*aktu&#xFFFD; (*aktu&#xFFFD; (*aktu&#xFFFD; (*aktu&#xFFFD; (*aktu&#xFFFD; (*aktu&#xFFFD; (*aktu&#xFFFD; (*aktu&#xFFFD; (*aktu&#xFFFD; (*aktu&#xFFFD; (*aktu&#xFFFD; (*aktu&#xFFFD; (*aktu&#xFFFD; (*aktu&#xFFFD; (*aktu&#xFFFD; (*aktu&#xFFFD; (*aktu&#xFFFD; (*aktu&#xFFFD; (*aktu&#xFFFD; (*aktu&#xFFFD; (*aktu&#xFFFD; (*aktu&#xFFFD; (*aktu&#xFFFD; (*aktu&#xFFFD; (*aktu&#xFFFD; (*aktu&#xFFFD; (*aktu&#xFFFD; (*aktu&#xFFFD; (*aktu&#xFFFD; (*aktu&#xFFFD; (*aktu&#xFFFD; (*aktu&#xFFFD; (*aktu&#xFFFD; (*aktu&#xFFFD; (*aktu&#xFFFD; (*aktu&#xFFFD; (*aktu&#xFFFD; (*aktu&#xFFFD; (*aktu&#xFFFD; (*aktu&#xFFFD; (*aktu&#xFFFD; (*aktu&#xFFFD; (*aktu&#xFFFD; (*aktu&#xFFFD; (*aktu&#xFFFD; (*aktu&#xFFFD; (*aktu&#xFFFD; (*aktu&#xFFFD; (*aktu&#xFFFD; (*aktu&#xFFFD; (*aktu&#xFFFD; (*aktu&#xFFFD; (*aktu&#xFFFD; (*aktu&#xFFFD; (*aktu&#xFFFD; (*aktu&#xFFFD; (*aktu&#xFFFD; (*aktu&#xFFFD; (*aktu&#xFFFD; (*aktu&#xFFFD; (*aktu&#xFFFD; (*aktu&#xFFFD; (*aktu&#xFFFD; (*aktu&#xFFFD; (*aktu&#xFFFD; (*aktu&#xFFFD; (*aktu&#xFFFD; (*aktu&#xFFFD; (*aktu&#xFFFD; (*aktu&#xFFFD; (*aktu&#xFFFD; (*aktu&#xFFFD; (*aktu&#xFFFD; (*aktu&#xFFFD; (*aktu&#xFFFD; (*aktu&#xFFFD; (*aktu&#xFFFD; (*aktu&#xFFFD; (*aktu&#xFFFD; (*aktu&#xFFFD; (*aktu&#xFFFD; (*aktu&#xFFFD; (*aktu&#xFFFD; (*aktu&#xFFFD; (*aktu&#xFFFD; (*aktu&#xFFFD; (*aktu&#xFFFD; (*aktu&#xFFFD; (*aktu&#xFFFD; (*aktu&#xFFFD; (*aktu&#xFFFD; (*aktu&#xFFFD; (*aktu&#xFFFD; (*aktu&#xFFFD; (*aktu&#xFFFD; (*aktu&#xFFFD; (*aktu&#xFFFD; (*aktu&#xFFFD; (*aktu&#xFFFD; (*aktu&#xFFFD; (*aktu&#xFFFD; (*aktu&#xFFFD; (*aktu&#xFFFD; (*aktu&#xFFFD; (*aktu&#xFFFD; (*aktu&#xFFFD; (*aktu&#xFFFD; (*aktu&#xFFFD; (*aktu&#xFFFD; (*aktu&#xFFFD; (*aktu&#xFFFD; (*aktu&#xFFFD; (*aktu&#xFFFD; (*aktu&#xFFFD; (*aktu&#xFFFD; (*aktu&#xFFFD; (*aktu&#xFFFD; (*aktu&#xFFFD; (*aktu&#xFFFD; (*aktu&#xFFFD; (*aktu&#xFFFD; (*aktu&#xFFFD; (*aktu&#xFFFD; (*aktu&#xFFFD; (*aktu&#xFFFD; (*aktu&#xFFFD; (*aktu&#xFFFD; (*aktu&#xFFFD; (*aktu&#xFFFD; (*aktu&#xFFFD; (*aktu&#xFFFD; (*aktu&#xFFFD; (*aktu&#xFFFD; (*aktu&#xFFFD; (*aktu&#xFFFD; (*aktu&#xFFFD; (*aktu&#xFFFD; (*aktu&#xFFFD; (*aktu&#xFFFD; (*aktu&#xFFFD; (*aktu&#xFFFD; (*aktu&#xFFFD; (*aktu&#xFFFD; (*aktu&#xFFFD; (*aktu&#xFFFD; (*aktu&#xFFFD; (*aktu&#xFFFD; (*aktu&#xFFFD; (*aktu&#xFFFD; (*aktu&#xFFFD; (*aktu&#xFFFD; (*aktu&#xFFFD; (*aktu&#xFFFD; (*aktu&#xFFFD; (*aktu&#xFFFD; (*aktu&#xFFFD; (*aktu&#xFFFD; (*aktu&#xFFFD; (*aktu&#xFFFD; (*aktu&#xFFFD; (*aktu&#xFFFD; (*aktu&#xFFFD; (*aktu&#xFFFD; (*aktu&#xFFFD; (*aktu&#xFFFD; (*aktu&#xFFFD; (*aktu&#xFFFD; (*aktu&#xFFFD; (*aktu&#xFFFD; (*aktu&#xFFFD; (*aktu&#xFFFD; (*aktu&#xFFFD; (*aktu&#xFFFD; (*aktu&#xFFFD; (*aktu&#xFFFD; (*aktu&#xFFFD; (*aktu&#xFFFD; (*aktu&#xFFFD; (*aktu&#xFFFD; (*aktu&#xFFFD; (*aktu&#xFFFD; (*aktu&#xFFFD; (*aktu&#xFFFD; (*aktu&#xFFFD; (*aktu&#xFFFD; (*aktu&#xFFFD; (*aktu&#xFFFD; (*aktu&#xFFFD; (*aktu&#xFFFD; (*aktu&#xFFFD; (*aktu&#xFFFD; (*aktu&#xFFFD; (*aktu&#xFFFD; (*aktu&#xFFFD; (*aktu&#xFFFD; (*aktu&#xFFFD; (*aktu&#xFFFD; (*aktu&#xFFFD; (*aktu&#xFFFD; (*aktu&#xFFFD; (*aktu&#xFFFD; (*aktu&#xFFFD; (*aktu&#xFFFD; (*aktu&#xFFFD; (*aktu&#xFFFD; (*aktu&#xFFFD; (*aktu&#xFFFD; (*aktu&#xFFFD; (*aktu&#xFFFD; (*aktu&#xFFFD; (*aktu&#xFFFD; (*aktu&#xFFFD; (*aktu&#xFFFD; (*aktu&#xFFFD; (*aktu&#xFFFD; (*aktu&#xFFFD; (*aktu&#xFFFD; (*aktu&#xFFFD; (*aktu&#xFFFD; (*aktu&#xFFFD; (*aktu&#xFFFD; (*aktu&#xFFFD; (*aktu&#xFFFD; (*aktu&#xFFFD; (*aktu&#xFFFD; (*aktu&#xFFFD; (*aktu&#xFFFD; (*aktu&#xFFFD; (*aktu&#xFFFD; (*aktu&#xFFFD; (*aktu&#xFFFD; (*aktu&#xFFFD; (*aktu&#xFFFD; (*aktu&#xFFFD; (*aktu&#xFFFD; (*aktu&#xFFFD; (*aktu&#xFFFD; (*aktu&#xFFFD; (*aktu&#xFFFD; (*aktu&#xFFFD; (*aktu&#xFFFD; (*aktu&#xFFFD; (*aktu&#xFFFD; (*aktu&#xFFFD; (*aktu&#xFFFD; (*aktu&#xFFFD; (*aktu&#xFFFD; (*aktu&#xFFFD; (*aktu&#xFFFD; (*aktu&#xFFFD; (*aktu&#xFFFD; (*aktu&#xFFFD; (*aktu&#xFFFD; (*aktu&#xFFFD; (*aktu&#xFFFD; (*aktu&#xFFFD; (*aktu&#xFFFD; (*aktu&#xFFFD; (*aktu&#xFFFD; (*aktu&#xFFFD; (*aktu&#xFFFD; (*aktu&#xFFFD; (*aktu&#xFFFD; (*aktu&#xFFFD; (*aktu&#xFFFD; (*aktu&#xFFFD; (*aktu&#xFFFD; (*aktu&#xFFFD; (*aktu&#xFFFD; (*aktu&#xFFFD; (*aktu&#xFFFD; (*aktu&#xFFFD; (*aktu&#xFFFD; (*aktu&#xFFFD; (*aktu&#xFFFD; (*aktu&#xFFFD; (*aktu&#xFFFD; (*aktu&#xFFFD; (*aktu&#xFFFD; (*aktu&#xFFFD; (*aktu&#xFFFD; (*aktu&#xFFFD; (*aktu&#xFFFD; (*aktu&#xFFFD; (*aktu&#xFFFD; (*aktu&#xFFFD; (*aktu&#xFFFD; (*aktu&#xFFFD; (*aktu&#xFFFD; (*aktu&#xFFFD; (*aktu&#xFFFD; (*aktu&#xFFFD; (*aktu&#xFFFD; (*aktu&#xFFFD; (*aktu&#xFFFD; (*aktu&#xFFFD; (*aktu&#xFFFD; (*aktu&#xFFFD; (*aktu&#xFFFD; (*aktu&#xFFFD; (*aktu&#xFFFD; (*aktu&#xFFFD; (*aktu&#xFFFD; (*aktu&#xFFFD; (*aktu&#xFFFD; (*aktu&#xFFFD; (*aktu&#xFFFD; (*aktu&#xFFFD; (*aktu&#xFFFD; (*aktu&#xFFFD; (*aktu&#xFFFD; (*aktu&#xFFFD; (*aktu&#xFFFD; (*aktu&#xFFFD; (*aktu&#xFFFD; (*aktu&#xFFFD; (*aktu&#xFFFD; (*aktu&#xFFFD; (*aktu&#xFFFD; (*aktu&#xFFFD; (*aktu&#xFFFD; (*aktu&#xFFFD; (*aktu&#xFFFD; (*aktu&#xFFFD; (*aktu&#xFFFD; (*aktu&#xFFFD; (*aktu&#xFFFD; (*aktu&#xFFFD; (*aktu&#xFFFD; (*aktu&#xFFFD; (*aktu&#xFFFD; (*aktu&#xFFFD; (*aktu&#xFFFD; (*aktu&#xFFFD; (*aktu&#xFFFD; (*aktu&#xFFFD; (*aktu&#xFFFD; (*aktu&#xFFFD; (*aktu&#xFFFD; (*aktu&#xFFFD; (*aktu&#xFFFD; (*aktu&#xFFFD; (*aktu&#xFFFD; (*aktu&#xFFFD; (*aktu&#xFFFD; (*aktu&#xFFFD; (*aktu&#xFFFD; (*aktu&#xFFFD; (*aktu&#xFFFD; (*aktu&#xFFFD; (*aktu&#xFFFD; (*aktu&#xFFFD; (*aktu&#xFFFD; (*aktu&#xFFFD; (*aktu&#xFFFD; (*aktu&#xFFFD; (*aktu&#xFFFD; (*aktu&#xFFFD; (*aktu&#xFFFD; (*aktu&#xFFFD; (*aktu&#xFFFD; (*aktu&#xFFFD; (*aktu&#xFFFD; (*aktu&#xFFFD; (*aktu&#xFFFD; (*aktu&#xFFFD; (*aktu&#xFFFD; (*aktu&#xFFFD; (*aktu&#xFFFD; (*aktu&#xFFFD; (*aktu&#xFFFD; (*aktu&#xFFFD; (*aktu&#xFFFD; (*aktu&#xFFFD; (*aktu&#xFFFD; (*aktu&#xFFFD; (*aktu&#xFFFD; (*aktu&#xFFFD; (*aktu&#xFFFD; (*aktu&#xFFFD; (*aktu&#xFFFD; (*aktu&#xFFFD; (*aktu&#xFFFD; (*aktu&#xFFFD; (*aktu&#xFFFD; (*aktu&#xFFFD; (*aktu&#xFFFD; (*aktu&#xFFFD; (*aktu&#xFFFD; (*aktu&#xFFFD; (*aktu&#xFFFD; (*aktu&#xFFFD; (*aktu&#xFFFD; (*aktu&#xFFFD; (*aktu&#xFFFD; (*aktu&#xFFFD; (*aktu&#xFFFD; (*aktu&#xFFFD; (*aktu&#xFFFD; (*aktu&#xFFFD; (*aktu&#xFFFD; (*aktu&#xFFFD; (*aktu&#xFFFD; (*aktu&#xFFFD; (*aktu&#xFFFD; (*aktu&#xFFFD; (*aktu&#xFFFD; (*aktu&#xFFFD; (*aktu&#xFFFD; (*aktu&#xFFFD; (*aktu&#xFFFD; (*aktu&#xFFFD; (*aktu&#xFFFD; (*aktu&#xFFFD; (*aktu&#xFFFD; (*aktu&#xFFFD; (*aktu&#xFFFD; (*aktu&#xFFFD; (*aktu&#xFFFD; (*aktu&#xFFFD; (*aktu&#xFFFD; (*aktu&#xFFFD; (*aktu&#xFFFD; (*aktu&#xFFFD; (*aktu&#xFFFD; (*aktu&#xFFFD; (*aktu&#xFFFD; (*aktu&#xFFFD; (*aktu&#xFFFD; (*aktu&#xFFFD; (*aktu&#xFFFD; (*aktu&#xFFFD; (*aktu&#xFFFD; (*aktu&#xFFFD; (*aktu&#xFFFD; (*aktu&#xFFFD; (*aktu&#xFFFD; (*aktu&#xFFFD; (*aktu&#xFFFD; (*aktu&#xFFFD; (*aktu&#xFFFD; (*aktu&#xFFFD; (*aktu&#xFFFD; (*aktu&#xFFFD; (*aktu&#xFFFD; (*aktu&#xFFFD; (*aktu&#xFFFD; (*aktu&#xFFFD; (*aktu&#xFFFD; (*aktu&#xFFFD; (*aktu&#xFFFD; (*aktu&#xFFFD; (*aktu&#xFFFD; (*aktu&#xFFFD; (*aktu&#xFFFD; (*aktu&#xFFFD; (*aktu&#xFFFD; (*aktu&#xFFFD; (*aktu&#xFFFD; (*aktu&#xFFFD; (*aktu&#xFFFD; (*aktu&#xFFFD; (*aktu&#xFFFD; (*aktu&#xFFFD; (*aktu&#xFFFD; (*aktu&#xFFFD; (*aktu&#xFFFD; (*aktu&#xFFFD; (*aktu&#xFFFD; (*aktu&#xFFFD; (*aktu&#xFFFD; (*aktu&#xFFFD; (*aktu&#xFFFD; (*aktu&#xFFFD; (*aktu&#xFFFD; (*aktu&#xFFFD; (*aktu&#xFFFD; (*aktu&#xFFFD; (*aktu&#xFFFD; (*aktu&#xFFFD; (*aktu&#xFFFD; (*aktu&#xFFFD; (*aktu&#xFFFD; (*aktu&#xFFFD; (*aktu&#xFFFD; (*aktu&#xFFFD; (*aktu&#xFFFD; (*aktu&#xFFFD; (*aktu&#xFFFD; (*aktu&#xFFFD; (*aktu&#xFFFD; (*aktu&#xFFFD; (*aktu&#xFFFD; (*aktu&#xFFFD; (*aktu&#xFFFD; (*aktu&#xFFFD; (*aktu&#xFFFD; (*aktu&#xFFFD; (*aktu&#xFFFD; (*aktu&#xFFFD; (*aktu&#xFFFD; (*aktu&#xFFFD; (*aktu&#xFFFD; (*aktu&#xFFFD; (*aktu&#xFFFD; (*aktu&#xFFFD; (*aktu&#xFFFD; (*aktu&#xFFFD; (*aktu&#xFFFD; (*aktu&#xFFFD; (*aktu&#xFFFD; (*aktu&#xFFFD; (*aktu&#xFFFD; (*aktu&#xFFFD; (*aktu&#xFFFD; (*aktu&#xFFFD; (*aktu&#xFFFD; (*aktu&#xFFFD; (*aktu&#xFFFD; (*aktu&#xFFFD; (*aktu&#xFFFD; (*aktu&#xFFFD; (*aktu&#xFFFD; (*aktu&#xFFFD; (*aktu&#xFFFD; (*aktu&#xFFFD; (*aktu&#xFFFD; (*aktu&#xFFFD; (*aktu&#xFFFD; (*aktu&#xFFFD; (*aktu&#xFFFD; (*aktu&#xFFFD; (*aktu&#xFFFD; (*aktu&#xFFFD; (*aktu&#xFFFD; (*aktu&#xFFFD; (*aktu&#xFFFD; (*aktu&#xFFFD; (*aktu&#xFFFD; (*aktu&#xFFFD; (*aktu&#xFFFD; (*aktu&#xFFFD; (*aktu&#xFFFD; (*aktu&#xFFFD; (*aktu&#xFFFD; (*aktu&#xFFFD; (*aktu&#xFFFD; (*aktu&#xFFFD; (*aktu&#xFFFD; (*aktu&#xFFFD; (*aktu&#xFFFD; (*aktu&#xFFFD; (*aktu&#xFFFD; (*aktu&#xFFFD; (*aktu&#xFFFD; (*aktu&#xFFFD; (*aktu&#xFFFD; (*aktu&#xFFFD; (*aktu&#xFFFD; (*aktu&#xFFFD; (*aktu&#xFFFD; (*aktu&#xFFFD; (*aktu&#xFFFD; (*aktu&#xFFFD; (*aktu&#xFFFD; (*aktu&#xFFFD; (*aktu&#xFFFD; (*aktu&#xFFFD; (*aktu&#xFFFD; (*aktu&#xFFFD; (*aktu&#xFFFD; (*aktu&#xFFFD; (*aktu&#xFFFD; (*aktu&#xFFFD; (*aktu&#xFFFD; (*aktu&#xFFFD; (*aktu&#xFFFD; (*aktu&#xFFFD; (*aktu&#xFFFD; (*aktu&#xFFFD; (*aktu&#xFFFD; (*aktu&#xFFFD; (*aktu&#xFFFD; (*aktu&#xFFFD; (*aktu&#xFFFD; (*aktu&#xFFFD; (*aktu&#xFFFD; (*aktu&#xFFFD; (*aktu&#xFFFD; (*aktu&#xFFFD; (*aktu&#xFFFD; (*aktu&#xFFFD; (*aktu&#xFFFD; (*aktu&#xFFFD; (*aktu&#xFFFD; (*aktu&#xFFFD; (*aktu&#xFFFD; (*aktu&#xFFFD; (*aktu&#xFFFD; (*aktu&#xFFFD; (*aktu&#xFFFD; (*aktu&#xFFFD; (*aktu&#xFFFD; (*aktu&#xFFFD; (*aktu&#xFFFD; (*aktu&#xFFFD; (*aktu&#xFFFD; (*aktu&#xFFFD; (*aktu&#xFFFD; (*aktu&#xFFFD; (*aktu&#xFFFD; (*aktu&#xFFFD; (*aktu&#xFFFD; (*aktu&#xFFFD; (*aktu&#xFFFD; (*aktu&#xFFFD; (*aktu&#xFFFD; (*aktu&#xFFFD; (*aktu&#xFFFD; (*aktu&#xFFFD; (*aktu&#xFFFD; (*aktu&#xFFFD; (*aktu&#xFFFD; (*aktu&#xFFFD; (*aktu&#xFFFD; (*aktu&#xFFFD; (*aktu&#xFFFD; (*aktu&#xFFFD; (*aktu&#xFFFD; (*aktu&#xFFFD; (*aktu&#xFFFD; (*aktu&#xFFFD; (*aktu&#xFFFD; (*aktu&#xFFFD; (*aktu&#xFFFD; (*aktu&#xFFFD; (*aktu&#xFFFD; (*aktu&#xFFFD; (*aktu&#xFFFD; (*aktu&#xFFFD; (*aktu&#xFFFD; (*aktu&#xFFFD; (*aktu&#xFFFD; (*aktu&#xFFFD; (*aktu&#xFFFD; (*aktu&#xFFFD; (*aktu&#xFFFD; (*aktu&#xFFFD; (*aktu&#xFFFD; (*aktu&#xFFFD; (*aktu&#xFFFD; (*aktu&#xFFFD; (*aktu&#xFFFD; (*aktu&#xFFFD; (*aktu&#xFFFD; (*aktu&#xFFFD; (*aktu&#xFFFD; (*aktu&#xFFFD; (*aktu&#xFFFD; (*aktu&#xFFFD; (*aktu&#xFFFD; (*aktu&#xFFFD; (*aktu&#xFFFD; (*aktu&#xFFFD; (*aktu&#xFFFD; (*aktu&#xFFFD; (*aktu&#xFFFD; (*aktu&#xFFFD; (*aktu&#xFFFD; (*aktu&#xFFFD; (*aktu&#xFFFD; (*aktu&#xFFFD; (*aktu&#xFFFD; (*aktu&#xFFFD; (*aktu&#xFFFD; (*aktu&#xFFFD; (*aktu&#xFFFD; (*aktu&#xFFFD; (*aktu&#xFFFD; (*aktu&#xFFFD; (*aktu&#xFFFD; (*aktu&#xFFFD; (*aktu&#xFFFD; (*aktu&#xFFFD; (*aktu&#xFFFD; (*aktu&#xFFFD; (*aktu&#xFFFD; (*aktu&#xFFFD; (*aktu&#xFFFD; (*aktu&#xFFFD; (*aktu&#xFFFD; (*aktu&#xFFFD; (*aktu&#xFFFD; (*aktu&#xFFFD; (*aktu&#xFFFD; (*aktu&#xFFFD; (*aktu&#xFFFD; (*aktu&#xFFFD; (*aktu&#xFFFD; (*aktu&#xFFFD; (*aktu&#xFFFD; (*aktu&#xFFFD; (*aktu&#xFFFD; (*aktu&#xFFFD; (*aktu&#xFFFD; (*aktu&#xFFFD; (*aktu&#xFFFD; (*aktu&#xFFFD; (*aktu&#xFFFD; (*aktu&#xFFFD; (*aktu&#xFFFD; (*aktu&#xFFFD; (*aktu&#xFFFD; (*aktu&#xFFFD; (*aktu&#xFFFD; (*aktu&#xFFFD; (*aktu&#xFFFD; (*aktu&#xFFFD; (*aktu&#xFFFD; (*aktu&#xFFFD; (*aktu&#xFFFD; (*aktu&#xFFFD; (*aktu&#xFFFD; (*aktu&#xFFFD; (*aktu&#xFFFD; (*aktu&#xFFFD; (*aktu&#xFFFD; (*aktu&#xFFFD; (*aktu&#xFFFD; (*aktu&#xFFFD; (*aktu&#xFFFD; (*aktu&#xFFFD; (*aktu&#xFFFD; (*aktu&#xFFFD; (*aktu&#xFFFD; (*aktu&#xFFFD; (*aktu&#xFFFD; (*aktu&#xFFFD; (*aktu&#xFFFD; (*aktu&#xFFFD; (*aktu&#xFFFD; (*aktu&#xFFFD; (*aktu&#xFFFD; (*aktu&#xFFFD; (*aktu&#xFFFD; (*aktu&#xFFFD; (*aktu&#xFFFD; (*aktu&#xFFFD; (*aktu&#xFFFD; (*aktu&#xFFFD; (*aktu&#xFFFD; (*aktu&#xFFFD; (*aktu&#xFFFD; (*aktu&#xFFFD; (*aktu&#xFFFD; (*aktu&#xFFFD; (*aktu&#xFFFD; (*aktu&#xFFFD; (*aktu&#xFFFD; (*aktu&#xFFFD; (*aktu&#xFFFD; (*aktu&#xFFFD; (*aktu&#xFFFD; (*aktu&#xFFFD; (*aktu&#xFFFD; (*aktu&#xFFFD; (*aktu&#xFFFD; (*aktu&#xFFFD; (*aktu&#xFFFD; (*aktu&#xFFFD; (*aktu&#xFFFD; (*aktu&#xFFFD; (*aktu&#xFFFD; (*aktu&#xFFFD; (*aktu&#xFFFD; (*aktu&#xFFFD; (*aktu&#xFFFD; (*aktu&#xFFFD; (*aktu&#xFFFD; (*aktu&#xFFFD; (*aktu&#xFFFD; (*aktu&#xFFFD; (*aktu&#xFFFD; (*aktu&#xFFFD; (*aktu&#xFFFD; (*aktu&#xFFFD; (*aktu&#xFFFD; (*aktu&#xFFFD; (*aktu&#xFFFD; (*aktu&#xFFFD; (*aktu&#xFFFD; (*aktu&#xFFFD; (*aktu&#xFFFD; (*aktu&#xFFFD; (*aktu&#xFFFD; (*aktu&#xFFFD; (*aktu&#xFFFD; (*aktu&#xFFFD; (*aktu&#xFFFD; (*aktu&#xFFFD; (*aktu&#xFFFD; (*aktu&#xFFFD; (*aktu&#xFFFD; (*aktu&#xFFFD; (*aktu&#xFFFD; (*aktu&#xFFFD; (*aktu&#xFFFD; (*aktu&#xFFFD; (*aktu&#xFFFD; (*aktu&#xFFFD; (*aktu&#xFFFD; (*aktu&#xFFFD; (*aktu&#xFFFD; (*aktu&#xFFFD; (*aktu&#xFFFD; (*aktu&#xFFFD; (*aktu&#xFFFD; (*aktu&#xFFFD; (*aktu&#xFFFD; (*aktu&#xFFFD; (*aktu&#xFFFD; (*aktu&#xFFFD; (*aktu&#xFFFD; (*aktu&#xFFFD; (*aktu&#xFFFD; (*aktu&#xFFFD; (*aktu&#xFFFD; (*aktu&#xFFFD; (*aktu&#xFFFD; (*aktu&#xFFFD; (*aktu&#xFFFD; (*aktu&#xFFFD; (*aktu&#xFFFD; (*aktu&#xFFFD; (*aktu&#xFFFD; (*aktu&#xFFFD; (*aktu&#xFFFD; (*aktu&#xFFFD; (*aktu&#xFFFD; (*aktu&#xFFFD; (*aktu&#xFFFD; (*aktu&#xFFFD; (*aktu&#xFFFD; (*aktu&#xFFFD; (*aktu&#xFFFD; (*aktu&#xFFFD; (*aktu&#xFFFD; (*aktu&#xFFFD; (*aktu&#xFFFD; (*aktu&#xFFFD; (*aktu&#xFFFD; (*aktu&#xFFFD; (*aktu&#xFFFD; (*aktu&#xFFFD; (*aktu&#xFFFD; (*aktu&#xFFFD; (*aktu&#xFFFD; (*aktu&#xFFFD; (*aktu&#xFFFD; (*aktu&#xFFFD; (*aktu&#xFFFD; (*aktu&#xFFFD; (*aktu&#xFFFD; (*aktu&#xFFFD; (*aktu&#xFFFD; (*aktu&#xFFFD; (*aktu&#xFFFD; (*aktu&#xFFFD; (*aktu&#xFFFD; (*aktu&#xFFFD; (*aktu&#xFFFD; (*aktu&#xFFFD; (*aktu&#xFFFD; (*aktu&#xFFFD; (*aktu&#xFFFD; (*aktu&#xFFFD; (*aktu&#xFFFD; (*aktu&#xFFFD; (*aktu&#xFFFD; (*aktu&#xFFFD; (*aktu&#xFFFD; (*aktu&#xFFFD; (*aktu&#xFFFD; (*aktu&#xFFFD; (*aktu&#xFFFD; (*aktu&#xFFFD; (*aktu&#xFFFD; (*aktu&#xFFFD; (*aktu&#xFFFD; (*aktu&#xFFFD; (*aktu&#xFFFD; (*aktu&#xFFFD; (*aktu&#xFFFD; (*aktu&#xFFFD; (*aktu&#xFFFD; (*aktu&#xFFFD; (*aktu&#xFFFD; (*aktu&#xFFFD; (*aktu&#xFFFD; (*aktu&#xFFFD; (*aktu&#xFFFD; (*aktu&#xFFFD; (*aktu&#xFFFD; (*aktu&#xFFFD; (*aktu&#xFFFD; (*aktu&#xFFFD; (*aktu&#xFFFD; (*aktu&#xFFFD; (*aktu&#xFFFD; (*aktu&#xFFFD; (*aktu&#xFFFD; (*aktu&#xFFFD; (*aktu&#xFFFD; (*aktu&#xFFFD; (*aktu&#xFFFD; (*aktu&#xFFFD; (*aktu&#xFFFD; (*aktu&#xFFFD; (*aktu&#xFFFD; (*aktu&#xFFFD; (*aktu&#xFFFD; (*aktu&#xFFFD; (*aktu&#xFFFD; (*aktu&#xFFFD; (*aktu&#xFFFD; (*aktu&#xFFFD; (*aktu&#xFFFD; (*aktu&#xFFFD; (*aktu&#xFFFD; (*aktu&#xFFFD; (*aktu&#xFFFD; (*aktu&#xFFFD; (*aktu&#xFFFD; (*aktu&#xFFFD; (*aktu&#xFFFD; (*aktu&#xFFFD; (*aktu&#xFFFD; (*aktu&#xFFFD; (*aktu&#xFFFD; (*aktu&#xFFFD; (*aktu&#xFFFD; (*aktu&#xFFFD; (*aktu&#xFFFD; (*aktu&#xFFFD; (*aktu&#xFFFD; (*aktu&#xFFFD; (*aktu&#xFFFD; (*aktu&#xFFFD; (*aktu&#xFFFD; (*aktu&#xFFFD; (*aktu&#xFFFD; (*aktu&#xFFFD; (*aktu&#xFFFD; (*aktu&#xFFFD; (*aktu&#xFFFD; (*aktu&#xFFFD; (*aktu&#xFFFD; (*aktu&#xFFFD; (*aktu&#xFFFD; (*aktu&#xFFFD; (*aktu&#xFFFD; (*aktu&#xFFFD; (*aktu&#xFFFD; (*aktu&#xFFFD; (*aktu&#xFFFD; (*aktu&#xFFFD; (*aktu&#xFFFD; (*aktu&#xFFFD; (*aktu&#xFFFD; (*aktu&#xFFFD; (*aktu&#xFFFD; (*aktu&#xFFFD; (*aktu&#xFFFD; (*aktu&#xFFFD; (*aktu&#xFFFD; (*aktu&#xFFFD; (*aktu&#xFFFD; (*aktu&#xFFFD; (*aktu&#xFFFD; (*aktu&#xFFFD; (*aktu&#xFFFD; (*aktu&#xFFFD; (*aktu&#xFFFD; (*aktu&#xFFFD; (*aktu&#xFFFD; (*aktu&#xFFFD; (*aktu&#xFFFD; (*aktu&#xFFFD; (*aktu&#xFFFD; (*aktu&#xFFFD; (*aktu&#xFFFD; (*aktu&#xFFFD; (*aktu&#xFFFD; (*aktu&#xFFFD; (*aktu&#xFFFD; (*aktu&#xFFFD; (*aktu&#xFFFD; (*aktu&#xFFFD; (*aktu&#xFFFD; (*aktu&#xFFFD; (*aktu&#xFFFD; (*aktu&#xFFFD; (*aktu&#xFFFD; (*aktu&#xFFFD; (*aktu&#xFFFD; (*aktu&#xFFFD; (*aktu&#xFFFD; (*aktu&#xFFFD; (*aktu&#xFFFD; (*aktu&#xFFFD; (*aktu&#xFFFD; (*aktu&#xFFFD; (*aktu&#xFFFD; (*aktu&#xFFFD; (*aktu&#xFFFD; (*aktu&#xFFFD; (*aktu&#xFFFD; (*aktu&#xFFFD; (*aktu&#xFFFD; (*aktu&#xFFFD; (*aktu&#xFFFD; (*aktu&#xFFFD; (*aktu&#xFFFD; (*aktu&#xFFFD; (*aktu&#xFFFD; (*aktu&#xFFFD; (*aktu&#xFFFD; (*aktu&#xFFFD; (*aktu&#xFFFD; (*aktu&#xFFFD; (*aktu&#xFFFD; (*aktu&#xFFFD; (*aktu&#xFFFD; (*aktu&#xFFFD; (*aktu&#xFFFD; (*aktu&#xFFFD; (*aktu&#xFFFD; (*aktu&#xFFFD; (*aktu&#xFFFD; (*aktu&#xFFFD; (*aktu&#xFFFD; (*aktu&#xFFFD; (*aktu&#xFFFD; (*aktu&#xFFFD; (*aktu&#xFFFD; (*aktu&#xFFFD; (*aktu&#xFFFD; (*aktu&#xFFFD; (*aktu&#xFFFD; (*aktu&#xFFFD; (*aktu&#xFFFD; (*aktu&#xFFFD; (*aktu&#xFFFD; (*aktu&#xFFFD; (*aktu&#xFFFD; (*aktu&#xFFFD; (*aktu&#xFFFD; (*aktu&#xFFFD; (*aktu&#xFFFD; (*aktu&#xFFFD; (*aktu&#xFFFD; (*aktu&#xFFFD; (*aktu&#xFFFD; (*aktu&#xFFFD; (*aktu&#xFFFD; (*aktu&#xFFFD; (*aktu&#xFFFD; (*aktu&#xFFFD; (*aktu&#xFFFD; (*aktu&#xFFFD; (*aktu&#xFFFD; (*aktu&#xFFFD; (*aktu&#xFFFD; (*aktu&#xFFFD; (*aktu&#xFFFD; (*aktu&#xFFFD; (*aktu&#xFFFD; (*aktu&#xFFFD; (*aktu&#xFFFD; (*aktu&#xFFFD; (*aktu&#xFFFD; (*aktu&#xFFFD; (*aktu&#xFFFD; (*aktu&#xFFFD; (*aktu&#xFFFD; (*aktu&#xFFFD; (*aktu&#xFFFD; (*aktu&#xFFFD; (*aktu&#xFFFD; (*aktu&#xFFFD; (*aktu&#xFFFD; (*aktu&#xFFFD; (*aktu&#xFFFD; (*aktu&#xFFFD; (*aktu&#xFFFD; (*aktu&#xFFFD; (*aktu&#xFFFD; (*aktu&#xFFFD; (*aktu&#xFFFD; (*aktu&#xFFFD; (*aktu&#xFFFD; (*aktu&#xFFFD; (*aktu&#xFFFD; (*aktu&#xFFFD; (*aktu&#xFFFD; (*aktu&#xFFFD; (*aktu&#xFFFD; (*aktu&#xFFFD; (*aktu&#xFFFD; (*aktu&#xFFFD; (*aktu&#xFFFD; (*aktu&#xFFFD; (*aktu&#xFFFD; (*aktu&#xFFFD; (*aktu&#xFFFD; (*aktu&#xFFFD; (*aktu&#xFFFD; (*aktu&#xFFFD; (*aktu&#xFFFD; (*aktu&#xFFFD; (*aktu&#xFFFD; (*aktu&#xFFFD; (*aktu&#xFFFD; (*aktu&#xFFFD; (*aktu&#xFFFD; (*aktu&#xFFFD; (*aktu&#xFFFD; (*aktu&#xFFFD; (*aktu&#xFFFD; (*aktu&#xFFFD; (*aktu&#xFFFD; (*aktu&#xFFFD; (*aktu&#xFFFD; (*aktu&#xFFFD; (*aktu&#xFFFD; (*aktu&#xFFFD; (*aktu&#xFFFD; (*aktu&#xFFFD; (*aktu&#xFFFD; (*aktu&#xFFFD; (*aktu&#xFFFD; (*aktu&#xFFFD; (*aktu&#xFFFD; (*aktu&#xFFFD; (*aktu&#xFFFD; (*aktu&#xFFFD; (*aktu&#xFFFD; (*aktu&#xFFFD; (*aktu&#xFFFD; (*aktu&#xFFFD; (*aktu&#xFFFD; (*aktu&#xFFFD; (*aktu&#xFFFD; (*aktu&#xFFFD; (*aktu&#xFFFD; (*aktu&#xFFFD; (*aktu&#xFFFD; (*aktu&#xFFFD; (*aktu&#xFFFD; (*aktu&#xFFFD; (*aktu&#xFFFD; (*aktu&#xFFFD; (*aktu&#xFFFD; (*aktu&#xFFFD; (*aktu&#xFFFD; (*aktu&#xFFFD; (*aktu&#xFFFD; (*aktu&#xFFFD; (*aktu&#xFFFD; (*aktu&#xFFFD; (*aktu&#xFFFD; (*aktu&#xFFFD; (*aktu&#xFFFD; (*aktu&#xFFFD; (*aktu&#xFFFD; (*aktu&#xFFFD; (*aktu&#xFFFD; (*aktu&#xFFFD; (*aktu&#xFFFD; (*aktu&#xFFFD; (*aktu&#xFFFD; (*aktu&#xFFFD; (*aktu&#xFFFD; (*aktu&#xFFFD; (*aktu&#xFFFD; (*aktu&#xFFFD; (*aktu&#xFFFD; (*aktu&#xFFFD; (*aktu&#xFFFD; (*aktu&#xFFFD; (*aktu&#xFFFD; (*aktu&#xFFFD; (*aktu&#xFFFD; (*aktu&#xFFFD; (*aktu&#xFFFD; (*aktu&#xFFFD; (*aktu&#xFFFD; (*aktu&#xFFFD; (*aktu&#xFFFD; (*aktu&#xFFFD; (*aktu&#xFFFD; (*aktu&#xFFFD; (*aktu&#xFFFD; (*aktu&#xFFFD; (*aktu&#xFFFD; (*aktu&#xFFFD; (*aktu&#xFFFD; (*aktu&#xFFFD; (*aktu&#xFFFD; (*aktu&#xFFFD; (*aktu&#xFFFD; (*aktu&#xFFFD; (*aktu&#xFFFD; (*aktu&#xFFFD; (*aktu&#xFFFD; (*aktu&#xFFFD; (*aktu&#xFFFD; (*aktu&#xFFFD; (*aktu&#xFFFD; (*aktu&#xFFFD; (*aktu&#xFFFD; (*aktu&#xFFFD; (*aktu&#xFFFD; (*aktu&#xFFFD; (*aktu&#xFFFD; (*aktu&#xFFFD; (*aktu&#xFFFD; (*aktu&#xFFFD; (*aktu&#xFFFD; (*aktu&#xFFFD; (*aktu&#xFFFD; (*aktu&#xFFFD; (*aktu&#xFFFD; (*aktu&#xFFFD; (*aktu&#xFFFD; (*aktu&#xFFFD; (*aktu&#xFFFD; (*aktu&#xFFFD; (*aktu&#xFFFD; (*aktu&#xFFFD; (*aktu&#xFFFD; (*aktu&#xFFFD; (*aktu&#xFFFD; (*aktu&#xFFFD; (*aktu&#xFFFD; (*aktu&#xFFFD; (*aktu&#xFFFD; (*aktu&#xFFFD; (*aktu&#xFFFD; (*aktu&#xFFFD; (*aktu&#xFFFD; (*aktu&#xFFFD; (*aktu&#xFFFD; (*aktu&#xFFFD; (*aktu&#xFFFD; (*aktu&#xFFFD; (*aktu&#xFFFD; (*aktu&#xFFFD; (*aktu&#xFFFD; (*aktu&#xFFFD; (*aktu&#xFFFD; (*aktu&#xFFFD; (*aktu&#xFFFD; (*aktu&#xFFFD; (*aktu&#xFFFD; (*aktu&#xFFFD; (*aktu&#xFFFD; (*aktu&#xFFFD; (*aktu&#xFFFD; (*aktu&#xFFFD; (*aktu&#xFFFD; (*aktu&#xFFFD; (*aktu&#xFFFD; (*aktu&#xFFFD; (*aktu&#xFFFD; (*aktu&#xFFFD; (*aktu&#xFFFD; (*aktu&#xFFFD; (*aktu&#xFFFD; (*aktu&#xFFFD; (*aktu&#xFFFD; (*aktu&#xFFFD; (*aktu&#xFFFD; (*aktu&#xFFFD; (*aktu&#xFFFD; (*aktu&#xFFFD; (*aktu&#xFFFD; (*aktu&#xFFFD; (*aktu&#xFFFD; (*aktu&#xFFFD; (*aktu&#xFFFD; (*aktu&#xFFFD; (*aktu&#xFFFD; (*aktu&#xFFFD; (*aktu&#xFFFD; (*aktu&#xFFFD; (*aktu&#xFFFD; (*aktu&#xFFFD; (*aktu&#xFFFD; (*aktu&#xFFFD; (*aktu&#xFFFD; (*aktu&#xFFFD; (*aktu&#xFFFD; (*aktu&#xFFFD; (*aktu&#xFFFD; (*aktu&#xFFFD; (*aktu&#xFFFD; (*aktu&#xFFFD; (*aktu&#xFFFD; (*aktu&#xFFFD; (*aktu&#xFFFD; (*aktu&#xFFFD; (*aktu&#xFFFD; (*aktu&#xFFFD; (*aktu&#xFFFD; (*aktu&#xFFFD; (*aktu&#xFFFD; (*aktu&#xFFFD; (*aktu&#xFFFD; (*aktu&#xFFFD; (*aktu&#xFFFD; (*aktu&#xFFFD; (*aktu&#xFFFD; (*aktu&#xFFFD; (*aktu&#xFFFD; (*aktu&#xFFFD; (*aktu&#xFFFD; (*aktu&#xFFFD; (*aktu&#xFFFD; (*aktu&#xFFFD; (*aktu&#xFFFD; (*aktu&#xFFFD; (*aktu&#xFFFD; (*aktu&#xFFFD; (*aktu&#xFFFD; (*aktu&#xFFFD; (*aktu&#xFFFD; (*aktu&#xFFFD; (*aktu&#xFFFD; (*aktu&#xFFFD; (*aktu&#xFFFD; (*aktu&#xFFFD; (*aktu&#xFFFD; (*aktu&#xFFFD; (*aktu&#xFFFD; (*aktu&#xFFFD; (*aktu&#xFFFD; (*aktu&#xFFFD; (*aktu&#xFFFD; (*aktu&#xFFFD; (*aktu&#xFFFD; (*aktu&#xFFFD; (*aktu&#xFFFD; (*aktu&#xFFFD; (*aktu&#xFFFD; (*aktu&#xFFFD; (*aktu&#xFFFD; (*aktu&#xFFFD; (*aktu&#xFFFD; (*aktu&#xFFFD; (*aktu&#xFFFD; (*aktu&#xFFFD; (*aktu&#xFFFD; (*aktu&#xFFFD; (*aktu&#xFFFD; (*aktu&#xFFFD; (*aktu&#xFFFD; (*aktu&#xFFFD; (*aktu&#xFFFD; (*aktu&#xFFFD; (*aktu&#xFFFD; (*aktu&#xFFFD; (*aktu&#xFFFD; (*aktu&#xFFFD; (*aktu&#xFFFD; (*aktu&#xFFFD; (*aktu&#xFFFD; (*aktu&#xFFFD; (*aktu&#xFFFD; (*aktu&#xFFFD; (*aktu&#xFFFD; (*aktu&#xFFFD; (*aktu&#xFFFD; (*aktu&#xFFFD; (*aktu&#xFFFD; (*aktu&#xFFFD; (*aktu&#xFFFD; (*aktu&#xFFFD; (*aktu&#xFFFD; (*aktu&#xFFFD; (*aktu&#xFFFD; (*aktu&#xFFFD; (*aktu&#xFFFD; (*aktu&#xFFFD; (*aktu&#xFFFD; (*aktu&#xFFFD; (*aktu&#xFFFD; (*aktu&#xFFFD; (*aktu&#xFFFD; (*aktu&#xFFFD; (*aktu&#xFFFD; (*aktu&#xFFFD; (*aktu&#xFFFD; (*aktu&#xFFFD; (*aktu&#xFFFD; (*aktu&#xFFFD; (*aktu&#xFFFD; (*aktu&#xFFFD; (*aktu&#xFFFD; (*aktu&#xFFFD; (*aktu&#xFFFD; (*aktu&#xFFFD; (*aktu&#xFFFD; (*aktu&#xFFFD; (*aktu&#xFFFD; (*aktu&#xFFFD; (*aktu&#xFFFD; (*aktu&#xFFFD; (*aktu&#xFFFD; (*aktu&#xFFFD; (*aktu&#xFFFD; (*aktu&#xFFFD; (*aktu&#xFFFD; (*aktu&#xFFFD; (*aktu&#xFFFD; (*aktu&#xFFFD; (*aktu&#xFFFD; (*aktu&#xFFFD; (*aktu&#xFFFD; (*aktu&#xFFFD; (*aktu&#xFFFD; (*aktu&#xFFFD; (*aktu&#xFFFD; (*aktu&#xFFFD; (*aktu&#xFFFD; (*aktu&#xFFFD; (*aktu&#xFFFD; (*aktu&#xFFFD; (*aktu&#xFFFD; (*aktu&#xFFFD; (*aktu&#xFFFD; (*aktu&#xFFFD; (*aktu&#xFFFD; (*aktu&#xFFFD; (*aktu&#xFFFD; (*aktu&#xFFFD; (*aktu&#xFFFD; (*aktu&#xFFFD; (*aktu&#xFFFD; (*aktu&#xFFFD; (*aktu&#xFFFD; (*aktu&#xFFFD; (*aktu&#xFFFD; (*aktu&#xFFFD; (*aktu&#xFFFD; (*aktu&#xFFFD; (*aktu&#xFFFD; (*aktu&#xFFFD; (*aktu&#xFFFD; (*aktu&#xFFFD; (*aktu&#xFFFD; (*aktu&#xFFFD; (*aktu&#xFFFD; (*aktu&#xFFFD; (*aktu&#xFFFD; (*aktu&#xFFFD; (*aktu&#xFFFD; (*aktu&#xFFFD; (*aktu&#xFFFD; (*aktu&#xFFFD; (*aktu&#xFFFD; (*aktu&#xFFFD; (*aktu&#xFFFD; (*aktu&#xFFFD; (*aktu&#xFFFD; (*aktu&#xFFFD; (*aktu&#xFFFD; (*aktu&#xFFFD; (*aktu&#xFFFD; (*aktu&#xFFFD; (*aktu&#xFFFD; (*aktu&#xFFFD; (*aktu&#xFFFD; (*aktu&#xFFFD; (*aktu&#xFFFD; (*aktu&#xFFFD; (*aktu&#xFFFD; (*aktu&#xFFFD; (*aktu&#xFFFD; (*aktu&#xFFFD; (*aktu&#xFFFD; (*aktu&#xFFFD; (*aktu&#xFFFD; (*aktu&#xFFFD; (*aktu&#xFFFD; (*aktu&#xFFFD; (*aktu&#xFFFD; (*aktu&#xFFFD; (*aktu&#xFFFD; (*aktu&#xFFFD; (*aktu&#xFFFD; (*aktu&#xFFFD; (*aktu&#xFFFD; (*aktu&#xFFFD; (*aktu&#xFFFD; (*aktu&#xFFFD; (*aktu&#xFFFD; (*aktu&#xFFFD; (*aktu&#xFFFD; (*aktu&#xFFFD; (*aktu&#xFFFD; (*aktu&#xFFFD; (*aktu&#xFFFD; (*aktu&#xFFFD; (*aktu&#xFFFD; (*aktu&#xFFFD; (*aktu&#xFFFD; (*aktu&#xFFFD; (*aktu&#xFFFD; (*aktu&#xFFFD; (*aktu&#xFFFD; (*aktu&#xFFFD; (*aktu&#xFFFD; (*aktu&#xFFFD; (*aktu&#xFFFD; (*aktu&#xFFFD; (*aktu&#xFFFD; (*aktu&#xFFFD; (*aktu&#xFFFD; (*aktu&#xFFFD; (*aktu&#xFFFD; (*aktu&#xFFFD; (*aktu&#xFFFD; (*aktu&#xFFFD; (*aktu&#xFFFD; (*aktu&#xFFFD; (*aktu&#xFFFD; (*aktu&#xFFFD; (*aktu&#xFFFD; (*aktu&#xFFFD; (*aktu&#xFFFD; (*aktu&#xFFFD; (*aktu&#xFFFD; (*aktu&#xFFFD; (*aktu&#xFFFD; (*aktu&#xFFFD; (*aktu&#xFFFD; (*aktu&#xFFFD; (*aktu&#xFFFD; (*aktu&#xFFFD; (*aktu&#xFFFD; (*aktu&#xFFFD; (*aktu&#xFFFD; (*aktu&#xFFFD; (*aktu&#xFFFD; (*aktu&#xFFFD; (*aktu&#xFFFD; (*aktu&#xFFFD; (*aktu&#xFFFD; (*aktu&#xFFFD; (*aktu&#xFFFD; (*aktu&#xFFFD; (*aktu&#xFFFD; (*aktu&#xFFFD; (*aktu&#xFFFD; (*aktu&#xFFFD; (*aktu&#xFFFD; (*aktu&#xFFFD; (*aktu&#xFFFD; (*aktu&#xFFFD; (*aktu&#xFFFD; (*aktu&#xFFFD; (*aktu&#xFFFD; (*aktu&#xFFFD; (*aktu&#xFFFD; (*aktu&#xFFFD; (*aktu&#xFFFD; (*aktu&#xFFFD; (*aktu&#xFFFD; (*aktu&#xFFFD; (*aktu&#xFFFD; (*aktu&#xFFFD; (*aktu&#xFFFD; (*aktu&#xFFFD; (*aktu&#xFFFD; (*aktu&#xFFFD; (*aktu&#xFFFD; (*aktu&#xFFFD; (*aktu&#xFFFD; (*aktu&#xFFFD; (*aktu&#xFFFD; (*aktu&#xFFFD; (*aktu&#xFFFD; (*aktu&#xFFFD; (*aktu&#xFFFD; (*aktu&#xFFFD; (*aktu&#xFFFD; (*aktu&#xFFFD; (*aktu&#xFFFD; (*aktu&#xFFFD; (*aktu&#xFFFD; (*aktu&#xFFFD; (*aktu&#xFFFD; (*aktu&#xFFFD; (*aktu&#xFFFD; (*aktu&#xFFFD; (*aktu&#xFFFD; (*aktu&#xFFFD; (*aktu&#xFFFD; (*aktu&#xFFFD; (*aktu&#xFFFD; (*aktu&#xFFFD; (*aktu&#xFFFD; (*aktu&#xFFFD; (*aktu&#xFFFD; (*aktu&#xFFFD; (*aktu&#xFFFD; (*aktu&#xFFFD; (*aktu&#xFFFD; (*aktu&#xFFFD; (*aktu&#xFFFD; (*aktu&#xFFFD; (*aktu&#xFFFD; (*aktu&#xFFFD; (*aktu&#xFFFD; (*aktu&#xFFFD; (*aktu&#xFFFD; (*aktu&#xFFFD; (*aktu&#xFFFD; (*aktu&#xFFFD; (*aktu&#xFFFD; (*aktu&#xFFFD; (*aktu&#xFFFD; (*aktu&#xFFFD; (*aktu&#xFFFD; (*aktu&#xFFFD; (*aktu&#xFFFD; (*aktu&#xFFFD; (*aktu&#xFFFD; (*aktu&#xFFFD; (*aktu&#xFFFD; (*aktu&#xFFFD; (*aktu&#xFFFD; (*aktu&#xFFFD; (*aktu&#xFFFD; (*aktu&#xFFFD; (*aktu&#xFFFD; (*aktu&#xFFFD; (*aktu&#xFFFD; (*aktu&#xFFFD; (*aktu&#xFFFD; (*aktu&#xFFFD; (*aktu&#xFFFD; (*aktu&#xFFFD; (*aktu&#xFFFD; (*aktu&#xFFFD; (*aktu&#xFFFD; (*aktu&#xFFFD; (*aktu&#xFFFD; (*aktu&#xFFFD; (*aktu&#xFFFD; (*aktu&#xFFFD; (*aktu&#xFFFD; (*aktu&#xFFFD; (*aktu&#xFFFD; (*aktu&#xFFFD; (*aktu&#xFFFD; (*aktu&#xFFFD; (*aktu&#xFFFD; (*aktu&#xFFFD; (*aktu&#xFFFD; (*aktu&#xFFFD; (*aktu&#xFFFD; (*aktu&#xFFFD; (*aktu&#xFFFD; (*aktu&#xFFFD; (*aktu&#xFFFD; (*aktu&#xFFFD; (*aktu&#xFFFD; (*aktu&#xFFFD; (*aktu&#xFFFD; (*aktu&#xFFFD; (*aktu&#xFFFD; (*aktu&#xFFFD; (*aktu&#xFFFD; (*aktu&#xFFFD; (*aktu&#xFFFD; (*aktu&#xFFFD; (*aktu&#xFFFD; (*aktu&#xFFFD; (*aktu&#xFFFD; (*aktu&#xFFFD; (*aktu&#xFFFD; (*aktu&#xFFFD; (*aktu&#xFFFD; (*aktu&#xFFFD; (*aktu&#xFFFD; (*aktu&#xFFFD; (*aktu&#xFFFD; (*aktu&#xFFFD; (*aktu&#xFFFD; (*aktu&#xFFFD; (*aktu&#xFFFD; (*aktu&#xFFFD; (*aktu&#xFFFD; (*aktu&#xFFFD; (*aktu&#xFFFD; (*aktu&#xFFFD; (*aktu&#xFFFD; (*aktu&#xFFFD; (*aktu&#xFFFD; (*aktu&#xFFFD; (*aktu&#xFFFD; (*aktu&#xFFFD; (*aktu&#xFFFD; (*aktu&#xFFFD; (*aktu&#xFFFD; (*aktu&#xFFFD; (*aktu&#xFFFD; (*aktu&#xFFFD; (*aktu&#xFFFD; (*aktu&#xFFFD; (*aktu&#xFFFD; (*aktu&#xFFFD; (*aktu&#xFFFD; (*aktu&#xFFFD; (*aktu&#xFFFD; (*aktu&#xFFFD; (*aktu&#xFFFD; (*aktu&#xFFFD; (*aktu&#xFFFD; (*aktu&#xFFFD; (*aktu&#xFFFD; (*aktu&#xFFFD; (*aktu&#xFFFD; (*aktu&#xFFFD; (*aktu&#xFFFD; (*aktu&#xFFFD; (*aktu&#xFFFD; (*aktu&#xFFFD; (*aktu&#xFFFD; (*aktu&#xFFFD; (*aktu&#xFFFD; (*aktu&#xFFFD; (*aktu&#xFFFD; (*aktu&#xFFFD; (*aktu&#xFFFD; (*aktu&#xFFFD; (*aktu&#xFFFD; (*aktu&#xFFFD; (*aktu&#xFFFD; (*aktu&#xFFFD; (*aktu&#xFFFD; (*aktu&#xFFFD; (*aktu&#xFFFD; (*aktu&#xFFFD; (*aktu&#xFFFD; (*aktu&#xFFFD; (*aktu&#xFFFD; (*aktu&#xFFFD; (*aktu&#xFFFD; (*aktu&#xFFFD; (*aktu&#xFFFD; (*aktu&#xFFFD; (*aktu&#xFFFD; (*aktu&#xFFFD; (*aktu&#xFFFD; (*aktu&#xFFFD; (*aktu&#xFFFD; (*aktu&#xFFFD; (*aktu&#xFFFD; (*aktu&#xFFFD; (*aktu&#xFFFD; (*aktu&#xFFFD; (*aktu&#xFFFD; (*aktu&#xFFFD; (*aktu&#xFFFD; (*aktu&#xFFFD; (*aktu&#xFFFD; (*aktu&#xFFFD; (*aktu&#xFFFD; (*aktu&#xFFFD; (*aktu&#xFFFD; (*aktu&#xFFFD; (*aktu&#xFFFD; (*aktu&#xFFFD; (*aktu&#xFFFD; (*aktu&#xFFFD; (*aktu&#xFFFD; (*aktu&#xFFFD; (*aktu&#xFFFD; (*aktu&#xFFFD; (*aktu&#xFFFD; (*aktu&#xFFFD; (*aktu&#xFFFD; (*aktu&#xFFFD; (*aktu&#xFFFD; (*aktu&#xFFFD; (*aktu&#xFFFD; (*aktu&#xFFFD; (*aktu&#xFFFD; (*aktu&#xFFFD; (*aktu&#xFFFD; (*aktu&#xFFFD; (*aktu&#xFFFD; (*aktu&#xFFFD; (*aktu&#xFFFD; (*aktu&#xFFFD; (*aktu&#xFFFD; (*aktu&#xFFFD; (*aktu&#xFFFD; (*aktu&#xFFFD; (*aktu&#xFFFD; (*aktu&#xFFFD; (*aktu&#xFFFD; (*aktu&#xFFFD; (*aktu&#xFFFD; (*aktu&#xFFFD; (*aktu&#xFFFD; (*aktu&#xFFFD; (*aktu&#xFFFD; (*aktu&#xFFFD; (*aktu&#xFFFD; (*aktu&#xFFFD; (*aktu&#xFFFD; (*aktu&#xFFFD; (*aktu&#xFFFD; (*aktu&#xFFFD; (*aktu&#xFFFD; (*aktu&#xFFFD; (*aktu&#xFFFD; (*aktu&#xFFFD; (*aktu&#xFFFD; (*aktu&#xFFFD; (*aktu&#xFFFD; (*aktu&#xFFFD; (*aktu&#xFFFD; (*aktu&#xFFFD; (*aktu&#xFFFD; (*aktu&#xFFFD; (*aktu&#xFFFD; (*aktu&#xFFFD; (*aktu&#xFFFD; (*aktu&#xFFFD; (*aktu&#xFFFD; (*aktu&#xFFFD; (*aktu&#xFFFD; (*aktu&#xFFFD; (*aktu&#xFFFD; (*aktu&#xFFFD; (*aktu&#xFFFD; (*aktu&#xFFFD; (*aktu&#xFFFD; (*aktu&#xFFFD; (*aktu&#xFFFD; (*aktu&#xFFFD; (*aktu&#xFFFD; (*aktu&#xFFFD; (*aktu&#xFFFD; (*aktu&#xFFFD; (*aktu&#xFFFD; (*aktu&#xFFFD; (*aktu&#xFFFD; (*aktu&#xFFFD; (*aktu&#xFFFD; (*aktu&#xFFFD; (*aktu&#xFFFD; (*aktu&#xFFFD; (*aktu&#xFFFD; (*aktu&#xFFFD; (*aktu&#xFFFD; (*aktu&#xFFFD; (*aktu&#xFFFD; (*aktu&#xFFFD; (*aktu&#xFFFD; (*aktu&#xFFFD; (*aktu&#xFFFD; (*aktu&#xFFFD; (*aktu&#xFFFD; (*aktu&#xFFFD; (*aktu&#xFFFD; (*aktu&#xFFFD; (*aktu&#xFFFD; (*aktu&#xFFFD; (*aktu&#xFFFD; (*aktu&#xFFFD; (*aktu&#xFFFD; (*aktu&#xFFFD; (*aktu&#xFFFD; (*aktu&#xFFFD; (*aktu&#xFFFD; (*aktu&#xFFFD; (*aktu&#xFFFD; (*aktu&#xFFFD; (*aktu&#xFFFD; (*aktu&#xFFFD; (*aktu&#xFFFD; (*aktu&#xFFFD; (*aktu&#xFFFD; (*aktu&#xFFFD; (*aktu&#xFFFD; (*aktu&#xFFFD; (*aktu&#xFFFD; (*aktu&#xFFFD; (*aktu&#xFFFD; (*aktu&#xFFFD; (*aktu&#xFFFD; (*aktu&#xFFFD; (*aktu&#xFFFD; (*aktu&#xFFFD; (*aktu&#xFFFD; (*aktu&#xFFFD; (*aktu&#xFFFD; (*aktu&#xFFFD; (*aktu&#xFFFD; (*aktu&#xFFFD; (*aktu&#xFFFD; (*aktu&#xFFFD; (*aktu&#xFFFD; (*aktu&#xFFFD; (*aktu&#xFFFD; (*aktu&#xFFFD; (*aktu&#xFFFD; (*aktu&#xFFFD; (*aktu&#xFFFD; (*aktu&#xFFFD; (*aktu&#xFFFD; (*aktu&#xFFFD; (*aktu&#xFFFD; (*aktu&#xFFFD; (*aktu&#xFFFD; (*aktu&#xFFFD; (*aktu&#xFFFD; (*aktu&#xFFFD; (*aktu&#xFFFD; (*aktu&#xFFFD; (*aktu&#xFFFD; (*aktu&#xFFFD; (*aktu&#xFFFD; (*aktu&#xFFFD; (*aktu&#xFFFD; (*aktu&#xFFFD; (*aktu&#xFFFD; (*aktu&#xFFFD; (*aktu&#xFFFD; (*aktu&#xFFFD; (*aktu&#xFFFD; (*aktu&#xFFFD; (*aktu&#xFFFD; (*aktu&#xFFFD; (*aktu&#xFFFD; (*aktu&#xFFFD; (*aktu&#xFFFD; (*aktu&#xFFFD; (*aktu&#xFFFD; (*aktu&#xFFFD; (*aktu&#xFFFD; (*aktu&#xFFFD; (*aktu&#xFFFD; (*aktu&#xFFFD; (*aktu&#xFFFD; (*aktu&#xFFFD; (*aktu&#xFFFD; (*aktu&#xFFFD; (*aktu&#xFFFD; (*aktu&#xFFFD; (*aktu&#xFFFD; (*aktu&#xFFFD; (*aktu&#xFFFD; (*aktu&#xFFFD; (*aktu&#xFFFD; (*aktu&#xFFFD; (*aktu&#xFFFD; (*aktu&#xFFFD; (*aktu&#xFFFD; (*aktu&#xFFFD; (*aktu&#xFFFD; (*aktu&#xFFFD; (*aktu&#xFFFD; (*aktu&#xFFFD; (*aktu&#xFFFD; (*aktu&#xFFFD; (*aktu&#xFFFD; (*aktu&#xFFFD; (*aktu&#xFFFD; (*aktu&#xFFFD; (*aktu&#xFFFD; (*aktu&#xFFFD; (*aktu&#xFFFD; (*aktu&#xFFFD; (*aktu&#xFFFD; (*aktu&#xFFFD; (*aktu&#xFFFD; (*aktu&#xFFFD; (*aktu&#xFFFD; (*aktu&#xFFFD; (*aktu&#xFFFD; (*aktu&#xFFFD; (*aktu&#xFFFD; (*aktu&#xFFFD; (*aktu&#xFFFD; (*aktu&#xFFFD; (*aktu&#xFFFD; (*aktu&#xFFFD; (*aktu&#xFFFD; (*aktu&#xFFFD; (*aktu&#xFFFD; (*aktu&#xFFFD; (*aktu&#xFFFD; (*aktu&#xFFFD; (*aktu&#xFFFD; (*aktu&#xFFFD; (*aktu&#xFFFD; (*aktu&#xFFFD; (*aktu&#xFFFD; (*aktu&#xFFFD; (*aktu&#xFFFD; (*aktu&#xFFFD; (*aktu&#xFFFD; (*aktu&#xFFFD; (*aktu&#xFFFD; (*aktu&#xFFFD; (*aktu&#xFFFD; (*aktu&#xFFFD; (*aktu&#xFFFD; (*aktu&#xFFFD; (*aktu&#xFFFD; (*aktu&#xFFFD; (*aktu&#xFFFD; (*aktu&#xFFFD; (*aktu&#xFFFD; (*aktu&#xFFFD; (*aktu&#xFFFD; (*aktu&#xFFFD; (*aktu&#xFFFD; (*aktu&#xFFFD; (*aktu&#xFFFD; (*aktu&#xFFFD; (*aktu&#xFFFD; (*aktu&#xFFFD; (*aktu&#xFFFD; (*aktu&#xFFFD; (*aktu&#xFFFD; (*aktu&#xFFFD; (*aktu&#xFFFD; (*aktu&#xFFFD; (*aktu&#xFFFD; (*aktu&#xFFFD; (*aktu&#xFFFD; (*aktu&#xFFFD; (*aktu&#xFFFD; (*aktu&#xFFFD; (*aktu&#xFFFD; (*aktu&#xFFFD; (*aktu&#xFFFD; (*aktu&#xFFFD; (*aktu&#xFFFD; (*aktu&#xFFFD; (*aktu&#xFFFD; (*aktu&#xFFFD; (*aktu&#xFFFD; (*aktu&#xFFFD; (*aktu&#xFFFD; (*aktu&#xFFFD; (*aktu&#xFFFD; (*aktu&#xFFFD; (*aktu&#xFFFD; (*aktu&#xFFFD; (*aktu&#xFFFD; (*aktu&#xFFFD; (*aktu&#xFFFD; (*aktu&#xFFFD; (*aktu&#xFFFD; (*aktu&#xFFFD; (*aktu&#xFFFD; (*aktu&#xFFFD; (*aktu&#xFFFD; (*aktu&#xFFFD; (*aktu&#xFFFD; (*aktu&#xFFFD; (*aktu&#xFFFD; (*aktu&#xFFFD; (*aktu&#xFFFD; (*aktu&#xFFFD; (*aktu&#xFFFD; (*aktu&#xFFFD; (*aktu&#xFFFD; (*aktu&#xFFFD; (*aktu&#xFFFD; (*aktu&#xFFFD; (*aktu&#xFFFD; (*aktu&#xFFFD; (*aktu&#xFFFD; (*aktu&#xFFFD; (*aktu&#xFFFD; (*aktu&#xFFFD; (*aktu&#xFFFD; (*aktu&#xFFFD; (*aktu&#xFFFD; (*aktu&#xFFFD; (*aktu&#xFFFD; (*aktu&#xFFFD; (*aktu&#xFFFD; (*aktu&#xFFFD; (*aktu&#xFFFD; (*aktu&#xFFFD; (*aktu&#xFFFD; (*aktu&#xFFFD; (*aktu&#xFFFD; (*aktu&#xFFFD; (*aktu&#xFFFD; (*aktu&#xFFFD; (*aktu&#xFFFD; (*aktu&#xFFFD; (*aktu&#xFFFD; (*aktu&#xFFFD; (*aktu&#xFFFD; (*aktu&#xFFFD; (*aktu&#xFFFD; (*aktu&#xFFFD; (*aktu&#xFFFD; (*aktu&#xFFFD; (*aktu&#xFFFD; (*aktu&#xFFFD; (*aktu&#xFFFD; (*aktu&#xFFFD; (*aktu&#xFFFD; (*aktu&#xFFFD; (*aktu&#xFFFD; (*aktu&#xFFFD; (*aktu&#xFFFD; (*aktu&#xFFFD; (*aktu&#xFFFD; (*aktu&#xFFFD; (*aktu&#xFFFD; (*aktu&#xFFFD; (*aktu&#xFFFD; (*aktu&#xFFFD; (*aktu&#xFFFD; (*aktu&#xFFFD; (*aktu&#xFFFD; (*aktu&#xFFFD; (*aktu&#xFFFD; (*aktu&#xFFFD; (*aktu&#xFFFD; (*aktu&#xFFFD; (*aktu&#xFFFD; (*aktu&#xFFFD; (*aktu&#xFFFD; (*aktu&#xFFFD; (*aktu&#xFFFD; (*aktu&#xFFFD; (*aktu&#xFFFD; (*aktu&#xFFFD; (*aktu&#xFFFD; (*aktu&#xFFFD; (*aktu&#xFFFD; (*aktu&#xFFFD; (*aktu&#xFFFD; (*aktu&#xFFFD; (*aktu&#xFFFD; (*aktu&#xFFFD; (*aktu&#xFFFD; (*aktu&#xFFFD; (*aktu&#xFFFD; (*aktu&#xFFFD; (*aktu&#xFFFD; (*aktu&#xFFFD; (*aktu&#xFFFD; (*aktu&#xFFFD; (*aktu&#xFFFD; (*aktu&#xFFFD; (*aktu&#xFFFD; (*aktu&#xFFFD; (*aktu&#xFFFD; (*aktu&#xFFFD; (*aktu&#xFFFD; (*aktu&#xFFFD; (*aktu&#xFFFD; (*aktu&#xFFFD; (*aktu&#xFFFD; (*aktu&#xFFFD; (*aktu&#xFFFD; (*aktu&#xFFFD; (*aktu&#xFFFD; (*aktu&#xFFFD; (*aktu&#xFFFD; (*aktu&#xFFFD; (*aktu&#xFFFD; (*aktu&#xFFFD; (*aktu&#xFFFD; (*aktu&#xFFFD; (*aktu&#xFFFD; (*aktu&#xFFFD; (*aktu&#xFFFD; (*aktu&#xFFFD; (*aktu&#xFFFD; (*aktu&#xFFFD; (*aktu&#xFFFD; (*aktu&#xFFFD; (*aktu&#xFFFD; (*aktu&#xFFFD; (*aktu&#xFFFD; (*aktu&#xFFFD; (*aktu&#xFFFD; (*aktu&#xFFFD; (*aktu&#xFFFD; (*aktu&#xFFFD; (*aktu&#xFFFD; (*aktu&#xFFFD; (*aktu&#xFFFD; (*aktu&#xFFFD; (*aktu&#xFFFD; (*aktu&#xFFFD; (*aktu&#xFFFD; (*aktu&#xFFFD; (*aktu&#xFFFD; (*aktu&#xFFFD; (*aktu&#xFFFD; (*aktu&#xFFFD; (*aktu&#xFFFD; (*aktu&#xFFFD; (*aktu&#xFFFD; (*aktu&#xFFFD; (*aktu&#xFFFD; (*aktu&#xFFFD; (*aktu&#xFFFD; (*aktu&#xFFFD; (*aktu&#xFFFD; (*aktu&#xFFFD; (*aktu&#xFFFD; (*aktu&#xFFFD; (*aktu&#xFFFD; (*aktu&#xFFFD; (*aktu&#xFFFD; (*aktu&#xFFFD; (*aktu&#xFFFD; (*aktu&#xFFFD; (*aktu&#xFFFD; (*aktu&#xFFFD; (*aktu&#xFFFD; (*aktu&#xFFFD; (*aktu&#xFFFD; (*aktu&#xFFFD; (*aktu&#xFFFD; (*aktu&#xFFFD; (*aktu&#xFFFD; (*aktu&#xFFFD; (*aktu&#xFFFD; (*aktu&#xFFFD; (*aktu&#xFFFD; (*aktu&#xFFFD; (*aktu&#xFFFD; (*aktu&#xFFFD; (*aktu&#xFFFD; (*aktu&#xFFFD; (*aktu&#xFFFD; (*aktu&#xFFFD; (*aktu&#xFFFD; (*aktu&#xFFFD; (*aktu&#xFFFD; (*aktu&#xFFFD; (*aktu&#xFFFD; (*aktu&#xFFFD; (*aktu&#xFFFD; (*aktu&#xFFFD; (*aktu&#xFFFD; (*aktu&#xFFFD; (*aktu&#xFFFD; (*aktu&#xFFFD; (*aktu&#xFFFD; (*aktu&#xFFFD; (*aktu&#xFFFD; (*aktu&#xFFFD; (*aktu&#xFFFD; (*aktu&#xFFFD; (*aktu&#xFFFD; (*aktu&#xFFFD; (*aktu&#xFFFD; (*aktu&#xFFFD; (*aktu&#xFFFD; (*aktu&#xFFFD; (*aktu&#xFFFD; (*aktu&#xFFFD; (*aktu&#xFFFD; (*aktu&#xFFFD; (*aktu&#xFFFD; (*aktu&#xFFFD; (*aktu&#xFFFD; (*aktu&#xFFFD; (*aktu&#xFFFD; (*aktu&#xFFFD; (*aktu&#xFFFD; (*aktu&#xFFFD; (*aktu&#xFFFD; (*aktu&#xFFFD; (*aktu&#xFFFD; (*aktu&#xFFFD; (*aktu&#xFFFD; (*aktu&#xFFFD; (*aktu&#xFFFD; (*aktu&#xFFFD; (*aktu&#xFFFD; (*aktu&#xFFFD; (*aktu&#xFFFD; (*aktu&#xFFFD; (*aktu&#xFFFD; (*aktu&#xFFFD; (*aktu&#xFFFD; (*aktu&#xFFFD; (*aktu&#xFFFD; (*aktu&#xFFFD; (*aktu&#xFFFD; (*aktu&#xFFFD; (*aktu&#xFFFD; (*aktu&#xFFFD; (*aktu&#xFFFD; (*aktu&#xFFFD; (*aktu&#xFFFD; (*aktu&#xFFFD; (*aktu&#xFFFD; (*aktu&#xFFFD; (*aktu&#xFFFD; (*aktu&#xFFFD; (*aktu&#xFFFD; (*aktu&#xFFFD; (*aktu&#xFFFD; (*aktu&#xFFFD; (*aktu&#xFFFD; (*aktu&#xFFFD; (*aktu&#xFFFD; (*aktu&#xFFFD; (*aktu&#xFFFD; (*aktu&#xFFFD; (*aktu&#xFFFD; (*aktu&#xFFFD; (*aktu&#xFFFD; (*aktu&#xFFFD; (*aktu&#xFFFD; (*aktu&#xFFFD; (*aktu&#xFFFD; (*aktu&#xFFFD; (*aktu&#xFFFD; (*aktu&#xFFFD; (*aktu&#xFFFD; (*aktu&#xFFFD; (*aktu&#xFFFD; (*aktu&#xFFFD; (*aktu&#xFFFD; (*aktu&#xFFFD; (*aktu&#xFFFD; (*aktu&#xFFFD; (*aktu&#xFFFD; (*aktu&#xFFFD; (*aktu&#xFFFD; (*aktu&#xFFFD; (*aktu&#xFFFD; (*aktu&#xFFFD; (*aktu&#xFFFD; (*aktu&#xFFFD; (*aktu&#xFFFD; (*aktu&#xFFFD; (*aktu&#xFFFD; (*aktu&#xFFFD; (*aktu&#xFFFD; (*aktu&#xFFFD; (*aktu&#xFFFD; (*aktu&#xFFFD; (*aktu&#xFFFD; (*aktu&#xFFFD; (*aktu&#xFFFD; (*aktu&#xFFFD; (*aktu&#xFFFD; (*aktu&#xFFFD; (*aktu&#xFFFD; (*aktu&#xFFFD; (*aktu&#xFFFD; (*aktu&#xFFFD; (*aktu&#xFFFD; (*aktu&#xFFFD; (*aktu&#xFFFD; (*aktu&#xFFFD; (*aktu&#xFFFD; (*aktu&#xFFFD; (*aktu&#xFFFD; (*aktu&#xFFFD; (*aktu&#xFFFD; (*aktu&#xFFFD; (*aktu&#xFFFD; (*aktu&#xFFFD; (*aktu&#xFFFD; (*aktu&#xFFFD; (*aktu&#xFFFD; (*aktu&#xFFFD; (*aktu&#xFFFD; (*aktu&#xFFFD; (*aktu&#xFFFD; (*aktu&#xFFFD; (*aktu&#xFFFD; (*aktu&#xFFFD; (*aktu&#xFFFD; (*aktu&#xFFFD; (*aktu&#xFFFD; (*aktu&#xFFFD; (*aktu&#xFFFD; (*aktu&#xFFFD; (*aktu&#xFFFD; (*aktu&#xFFFD; (*aktu&#xFFFD; (*aktu&#xFFFD; (*aktu&#xFFFD; (*aktu&#xFFFD; (*aktu&#xFFFD; (*aktu&#xFFFD; (*aktu&#xFFFD; (*aktu&#xFFFD; (*aktu&#xFFFD; (*aktu&#xFFFD; (*aktu&#xFFFD; (*aktu&#xFFFD; (*aktu&#xFFFD; (*aktu&#xFFFD; (*aktu&#xFFFD; (*aktu&#xFFFD; (*aktu&#xFFFD; (*aktu&#xFFFD; (*aktu&#xFFFD; (*aktu&#xFFFD; (*aktu&#xFFFD; (*aktu&#xFFFD; (*aktu&#xFFFD; (*aktu&#xFFFD; (*aktu&#xFFFD; (*aktu&#xFFFD; (*aktu&#xFFFD; (*aktu&#xFFFD; (*aktu&#xFFFD; (*aktu&#xFFFD; (*aktu&#xFFFD; (*aktu&#xFFFD; (*aktu&#xFFFD; (*aktu&#xFFFD; (*aktu&#xFFFD; (*aktu&#xFFFD; (*aktu&#xFFFD; (*aktu&#xFFFD; (*aktu&#xFFFD; (*aktu&#xFFFD; (*aktu&#xFFFD; (*aktu&#xFFFD; (*aktu&#xFFFD; (*aktu&#xFFFD; (*aktu&#xFFFD; (*aktu&#xFFFD; (*aktu&#xFFFD; (*aktu&#xFFFD; (*aktu&#xFFFD; (*aktu&#xFFFD; (*aktu&#xFFFD; (*aktu&#xFFFD; (*aktu&#xFFFD; (*aktu&#xFFFD; (*aktu&#xFFFD; (*aktu&#xFFFD; (*aktu&#xFFFD; (*aktu&#xFFFD; (*aktu&#xFFFD; (*aktu&#xFFFD; (*aktu&#xFFFD; (*aktu&#xFFFD; (*aktu&#xFFFD; (*aktu&#xFFFD; (*aktu&#xFFFD; (*aktu&#xFFFD; (*aktu&#xFFFD; (*aktu&#xFFFD; (*aktu&#xFFFD; (*aktu&#xFFFD; (*aktu&#xFFFD; (*aktu&#xFFFD; (*aktu&#xFFFD; (*aktu&#xFFFD; (*aktu&#xFFFD; (*aktu&#xFFFD; (*aktu&#xFFFD; (*aktu&#xFFFD; (*aktu&#xFFFD; (*aktu&#xFFFD; (*aktu&#xFFFD; (*aktu&#xFFFD; (*aktu&#xFFFD; (*aktu&#xFFFD; (*aktu&#xFFFD; (*aktu&#xFFFD; (*aktu&#xFFFD; (*aktu&#xFFFD; (*aktu&#xFFFD; (*aktu&#xFFFD; (*aktu&#xFFFD; (*aktu&#xFFFD; (*aktu&#xFFFD; (*aktu&#xFFFD; (*aktu&#xFFFD; (*aktu&#xFFFD; (*aktu&#xFFFD; (*aktu&#xFFFD; (*aktu&#xFFFD; (*aktu&#xFFFD; (*aktu&#xFFFD; (*aktu&#xFFFD; (*aktu&#xFFFD; (*aktu&#xFFFD; (*aktu&#xFFFD; (*aktu&#xFFFD; (*aktu&#xFFFD; (*aktu&#xFFFD; (*aktu&#xFFFD; (*aktu&#xFFFD; (*aktu&#xFFFD; (*aktu&#xFFFD; (*aktu&#xFFFD; (*aktu&#xFFFD; (*aktu&#xFFFD; (*aktu&#xFFFD; (*aktu&#xFFFD; (*aktu&#xFFFD; (*aktu&#xFFFD; (*aktu&#xFFFD; (*aktu&#xFFFD; (*aktu&#xFFFD; (*aktu&#xFFFD; (*aktu&#xFFFD; (*aktu&#xFFFD; (*aktu&#xFFFD; (*aktu&#xFFFD; (*aktu&#xFFFD; (*aktu&#xFFFD; (*aktu&#xFFFD; (*aktu&#xFFFD; (*aktu&#xFFFD; (*aktu&#xFFFD; (*aktu&#xFFFD; (*aktu&#xFFFD; (*aktu&#xFFFD; (*aktu&#xFFFD; (*aktu&#xFFFD; (*aktu&#xFFFD; (*aktu&#xFFFD; (*aktu&#xFFFD; (*aktu&#xFFFD; (*aktu&#xFFFD; (*aktu&#xFFFD; (*aktu&#xFFFD; (*aktu&#xFFFD; (*aktu&#xFFFD; (*aktu&#xFFFD; (*aktu&#xFFFD; (*aktu&#xFFFD; (*aktu&#xFFFD; (*aktu&#xFFFD; (*aktu&#xFFFD; (*aktu&#xFFFD; (*aktu&#xFFFD; (*aktu&#xFFFD; (*aktu&#xFFFD; (*aktu&#xFFFD; (*aktu&#xFFFD; (*aktu&#xFFFD; (*aktu&#xFFFD; (*aktu&#xFFFD; (*aktu&#xFFFD; (*aktu&#xFFFD; (*aktu&#xFFFD; (*aktu&#xFFFD; (*aktu&#xFFFD; (*aktu&#xFFFD; (*aktu&#xFFFD; (*aktu&#xFFFD; (*aktu&#xFFFD; (*aktu&#xFFFD; (*aktu&#xFFFD; (*aktu&#xFFFD; (*aktu&#xFFFD; (*aktu&#xFFFD; (*aktu&#xFFFD; (*aktu&#xFFFD; (*aktu&#xFFFD; (*aktu&#xFFFD; (*aktu&#xFFFD; (*aktu&#xFFFD; (*aktu&#xFFFD; (*aktu&#xFFFD; (*aktu&#xFFFD; (*aktu&#xFFFD; (*aktu&#xFFFD; (*aktu&#xFFFD; (*aktu&#xFFFD; (*aktu&#xFFFD; (*aktu&#xFFFD; (*aktu&#xFFFD; (*aktu&#xFFFD; (*aktu&#xFFFD; (*aktu&#xFFFD; (*aktu&#xFFFD; (*aktu&#xFFFD; (*aktu&#xFFFD; (*aktu&#xFFFD; (*aktu&#xFFFD; (*aktu&#xFFFD; (*aktu&#xFFFD; (*aktu&#xFFFD; (*aktu&#xFFFD; (*aktu&#xFFFD; (*aktu&#xFFFD; (*aktu&#xFFFD; (*aktu&#xFFFD; (*aktu&#xFFFD; (*aktu&#xFFFD; (*aktu&#xFFFD; (*aktu&#xFFFD; (*aktu&#xFFFD; (*aktu&#xFFFD; (*aktu&#xFFFD; (*aktu&#xFFFD; (*aktu&#xFFFD; (*aktu&#xFFFD; (*aktu&#xFFFD; (*aktu&#xFFFD; (*aktu&#xFFFD; (*aktu&#xFFFD; (*aktu&#xFFFD; (*aktu&#xFFFD; (*aktu&#xFFFD; (*aktu&#xFFFD; (*aktu&#xFFFD; (*aktu&#xFFFD; (*aktu&#xFFFD; (*aktu&#xFFFD; (*aktu&#xFFFD; (*aktu&#xFFFD; (*aktu&#xFFFD; (*aktu&#xFFFD; (*aktu&#xFFFD; (*aktu&#xFFFD; (*aktu&#xFFFD; (*aktu&#xFFFD; (*aktu&#xFFFD; (*aktu&#xFFFD; (*aktu&#xFFFD; (*aktu&#xFFFD; (*aktu&#xFFFD; (*aktu&#xFFFD; (*aktu&#xFFFD; (*aktu&#xFFFD; (*aktu&#xFFFD; (*aktu&#xFFFD; (*aktu&#xFFFD; (*aktu&#xFFFD; (*aktu&#xFFFD; (*aktu&#xFFFD; (*aktu&#xFFFD; (*aktu&#xFFFD; (*aktu&#xFFFD; (*aktu&#xFFFD; (*aktu&#xFFFD; (*aktu&#xFFFD; (*aktu&#xFFFD; (*aktu&#xFFFD; (*aktu&#xFFFD; (*aktu&#xFFFD; (*aktu&#xFFFD; (*aktu&#xFFFD; (*aktu&#xFFFD; (*aktu&#xFFFD; (*aktu&#xFFFD; (*aktu&#xFFFD; (*aktu&#xFFFD; (*aktu&#xFFFD; (*aktu&#xFFFD; (*aktu&#xFFFD; (*aktu&#xFFFD; (*aktu&#xFFFD; (*aktu&#xFFFD; (*aktu&#xFFFD; (*aktu&#xFFFD; (*aktu&#xFFFD; (*aktu&#xFFFD; (*aktu&#xFFFD; (*aktu&#xFFFD; (*aktu&#xFFFD; (*aktu&#xFFFD; (*aktu&#xFFFD; (*aktu&#xFFFD; (*aktu&#xFFFD; (*aktu&#xFFFD; (*aktu&#xFFFD; (*aktu&#xFFFD; (*aktu&#xFFFD; (*aktu&#xFFFD; (*aktu&#xFFFD; (*aktu&#xFFFD; (*aktu&#xFFFD; (*aktu&#xFFFD; (*aktu&#xFFFD; (*aktu&#xFFFD; (*aktu&#xFFFD; (*aktu&#xFFFD; (*aktu&#xFFFD; (*aktu&#xFFFD; (*aktu&#xFFFD; (*aktu&#xFFFD; (*aktu&#xFFFD; (*aktu&#xFFFD; (*aktu&#xFFFD; (*aktu&#xFFFD; (*aktu&#xFFFD; (*aktu&#xFFFD; (*aktu&#xFFFD; (*aktu&#xFFFD; (*aktu&#xFFFD; (*aktu&#xFFFD; (*aktu&#xFFFD; (*aktu&#xFFFD; (*aktu&#xFFFD; (*aktu&#xFFFD; (*aktu&#xFFFD; (*aktu&#xFFFD; (*aktu&#xFFFD; (*aktu&#xFFFD; (*aktu&#xFFFD; (*aktu&#xFFFD; (*aktu&#xFFFD; (*aktu&#xFFFD; (*aktu&#xFFFD; (*aktu&#xFFFD; (*aktu&#xFFFD; (*aktu&#xFFFD; (*aktu&#xFFFD; (*aktu&#xFFFD; (*aktu&#xFFFD; (*aktu&#xFFFD; (*aktu&#xFFFD; (*aktu&#xFFFD; (*aktu&#xFFFD; (*aktu&#xFFFD; (*aktu&#xFFFD; (*aktu&#xFFFD; (*aktu&#xFFFD; (*aktu&#xFFFD; (*aktu&#xFFFD; (*aktu&#xFFFD; (*aktu&#xFFFD; (*aktu&#xFFFD; (*aktu&#xFFFD; (*aktu&#xFFFD; (*aktu&#xFFFD; (*aktu&#xFFFD; (*aktu&#xFFFD; (*aktu&#xFFFD; (*aktu&#xFFFD; (*aktu&#xFFFD; (*aktu&#xFFFD; (*aktu&#xFFFD; (*aktu&#xFFFD; (*aktu&#xFFFD; (*aktu&#xFFFD; (*aktu&#xFFFD; (*aktu&#xFFFD; (*aktu&#xFFFD; (*aktu&#xFFFD; (*aktu&#xFFFD; (*aktu&#xFFFD; (*aktu&#xFFFD; (*aktu&#xFFFD; (*aktu&#xFFFD; (*aktu&#xFFFD; (*aktu&#xFFFD; (*aktu&#xFFFD; (*aktu&#xFFFD; (*aktu&#xFFFD; (*aktu&#xFFFD; (*aktu&#xFFFD; (*aktu&#xFFFD; (*aktu&#xFFFD; (*aktu&#xFFFD; (*aktu&#xFFFD; (*aktu&#xFFFD; (*aktu&#xFFFD; (*aktu&#xFFFD; (*aktu&#xFFFD; (*aktu&#xFFFD; (*aktu&#xFFFD; (*aktu&#xFFFD; (*aktu&#xFFFD; (*aktu&#xFFFD; (*aktu&#xFFFD; (*aktu&#xFFFD; (*aktu&#xFFFD; (*aktu&#xFFFD; (*aktu&#xFFFD; (*aktu&#xFFFD; (*aktu&#xFFFD; (*aktu&#xFFFD; (*aktu&#xFFFD; (*aktu&#xFFFD; (*aktu&#xFFFD; (*aktu&#xFFFD; (*aktu&#xFFFD; (*aktu&#xFFFD; (*aktu&#xFFFD; (*aktu&#xFFFD; (*aktu&#xFFFD; (*aktu&#xFFFD; (*aktu&#xFFFD; (*aktu&#xFFFD; (*aktu&#xFFFD; (*aktu&#xFFFD; (*aktu&#xFFFD; (*aktu&#xFFFD; (*aktu&#xFFFD; (*aktu&#xFFFD; (*aktu&#xFFFD; (*aktu&#xFFFD; (*aktu&#xFFFD; (*aktu&#xFFFD; (*aktu&#xFFFD; (*aktu&#xFFFD; (*aktu&#xFFFD; (*aktu&#xFFFD; (*aktu&#xFFFD; (*aktu&#xFFFD; (*aktu&#xFFFD; (*aktu&#xFFFD; (*aktu&#xFFFD; (*aktu&#xFFFD; (*aktu&#xFFFD; (*aktu&#xFFFD; (*aktu&#xFFFD; (*aktu&#xFFFD; (*aktu&#xFFFD; (*aktu&#xFFFD; (*aktu&#xFFFD; (*aktu&#xFFFD; (*aktu&#xFFFD; (*aktu&#xFFFD; (*aktu&#xFFFD; (*aktu&#xFFFD; (*aktu&#xFFFD; (*aktu&#xFFFD; (*aktu&#xFFFD; (*aktu&#xFFFD; (*aktu&#xFFFD; (*aktu&#xFFFD; (*aktu&#xFFFD; (*aktu&#xFFFD; (*aktu&#xFFFD; (*aktu&#xFFFD; (*aktu&#xFFFD; (*aktu&#xFFFD; (*aktu&#xFFFD; (*aktu&#xFFFD; (*aktu&#xFFFD; (*aktu&#xFFFD; (*aktu&#xFFFD; (*aktu&#xFFFD; (*aktu&#xFFFD; (*aktu&#xFFFD; (*aktu&#xFFFD; (*aktu&#xFFFD; (*aktu&#xFFFD; (*aktu&#xFFFD; (*aktu&#xFFFD; (*aktu&#xFFFD; (*aktu&#xFFFD; (*aktu&#xFFFD; (*aktu&#xFFFD; (*aktu&#xFFFD; (*aktu&#xFFFD; (*aktu&#xFFFD; (*aktu&#xFFFD; (*aktu&#xFFFD; (*aktu&#xFFFD; (*aktu&#xFFFD; (*aktu&#xFFFD; (*aktu&#xFFFD; (*aktu&#xFFFD; (*aktu&#xFFFD; (*aktu&#xFFFD; (*aktu&#xFFFD; (*aktu&#xFFFD; (*aktu&#xFFFD; (*aktu&#xFFFD; (*aktu&#xFFFD; (*aktu&#xFFFD; (*aktu&#xFFFD; (*aktu&#xFFFD; (*aktu&#xFFFD; (*aktu&#xFFFD; (*aktu&#xFFFD; (*aktu&#xFFFD; (*aktu&#xFFFD; (*aktu&#xFFFD; (*aktu&#xFFFD; (*aktu&#xFFFD; (*aktu&#xFFFD; (*aktu&#xFFFD; (*aktu&#xFFFD; (*aktu&#xFFFD; (*aktu&#xFFFD; (*aktu&#xFFFD; (*aktu&#xFFFD; (*aktu&#xFFFD; (*aktu&#xFFFD; (*aktu&#xFFFD; (*aktu&#xFFFD; (*aktu&#xFFFD; (*aktu&#xFFFD; (*aktu&#xFFFD; (*aktu&#xFFFD; (*aktu&#xFFFD; (*aktu&#xFFFD; (*aktu&#xFFFD; (*aktu&#xFFFD; (*aktu&#xFFFD; (*aktu&#xFFFD; (*aktu&#xFFFD; (*aktu&#xFFFD; (*aktu&#xFFFD; (*aktu&#xFFFD; (*aktu&#xFFFD; (*aktu&#xFFFD; (*aktu&#xFFFD; (*aktu&#xFFFD; (*aktu&#xFFFD; (*aktu&#xFFFD; (*aktu&#xFFFD; (*aktu&#xFFFD; (*aktu&#xFFFD; (*aktu&#xFFFD; (*aktu&#xFFFD; (*aktu&#xFFFD; (*aktu&#xFFFD; (*aktu&#xFFFD; (*aktu&#xFFFD; (*aktu&#xFFFD; (*aktu&#xFFFD; (*aktu&#xFFFD; (*aktu&#xFFFD; (*aktu&#xFFFD; (*aktu&#xFFFD; (*aktu&#xFFFD; (*aktu&#xFFFD; (*aktu&#xFFFD; (*aktu&#xFFFD; (*aktu&#xFFFD; (*aktu&#xFFFD; (*aktu&#xFFFD; (*aktu&#xFFFD; (*aktu&#xFFFD; (*aktu&#xFFFD; (*aktu&#xFFFD; (*aktu&#xFFFD; (*aktu&#xFFFD; (*aktu&#xFFFD; (*aktu&#xFFFD; (*aktu&#xFFFD; (*aktu&#xFFFD; (*aktu&#xFFFD; (*aktu&#xFFFD; (*aktu&#xFFFD; (*aktu&#xFFFD; (*aktu&#xFFFD; (*aktu&#xFFFD; (*aktu&#xFFFD; (*aktu&#xFFFD; (*aktu&#xFFFD; (*aktu&#xFFFD; (*aktu&#xFFFD; (*aktu&#xFFFD; (*aktu&#xFFFD; (*aktu&#xFFFD; (*aktu&#xFFFD; (*aktu&#xFFFD; (*aktu&#xFFFD; (*aktu&#xFFFD; (*aktu&#xFFFD; (*aktu&#xFFFD; (*aktu&#xFFFD; (*aktu&#xFFFD; (*aktu&#xFFFD; (*aktu&#xFFFD; (*aktu&#xFFFD; (*aktu&#xFFFD; (*aktu&#xFFFD; (*aktu&#xFFFD; (*aktu&#xFFFD; (*aktu&#xFFFD; (*aktu&#xFFFD; (*aktu&#xFFFD; (*aktu&#xFFFD; (*aktu&#xFFFD; (*aktu&#xFFFD; (*aktu&#xFFFD; (*aktu&#xFFFD; (*aktu&#xFFFD; (*aktu&#xFFFD; (*aktu&#xFFFD; (*aktu&#xFFFD; (*aktu&#xFFFD; (*aktu&#xFFFD; (*aktu&#xFFFD; (*aktu&#xFFFD; (*aktu&#xFFFD; (*aktu&#xFFFD; (*aktu&#xFFFD; (*aktu&#xFFFD; (*aktu&#xFFFD; (*aktu&#xFFFD; (*aktu&#xFFFD; (*aktu&#xFFFD; (*aktu&#xFFFD; (*aktu&#xFFFD; (*aktu&#xFFFD; (*aktu&#xFFFD; (*aktu&#xFFFD; (*aktu&#xFFFD; (*aktu&#xFFFD; (*aktu&#xFFFD; (*aktu&#xFFFD; (*aktu&#xFFFD; (*aktu&#xFFFD; (*aktu&#xFFFD; (*aktu&#xFFFD; (*aktu&#xFFFD; (*aktu&#xFFFD; (*aktu&#xFFFD; (*aktu&#xFFFD; (*aktu&#xFFFD; (*aktu&#xFFFD; (*aktu&#xFFFD; (*aktu&#xFFFD; (*aktu&#xFFFD; (*aktu&#xFFFD; (*aktu&#xFFFD; (*aktu&#xFFFD; (*aktu&#xFFFD; (*aktu&#xFFFD; (*aktu&#xFFFD; (*aktu&#xFFFD; (*aktu&#xFFFD; (*aktu&#xFFFD; (*aktu&#xFFFD; (*aktu&#xFFFD; (*aktu&#xFFFD; (*aktu&#xFFFD; (*aktu&#xFFFD; (*aktu&#xFFFD; (*aktu&#xFFFD; (*aktu&#xFFFD; (*aktu&#xFFFD; (*aktu&#xFFFD; (*aktu&#xFFFD; (*aktu&#xFFFD; (*aktu&#xFFFD; (*aktu&#xFFFD; (*aktu&#xFFFD; (*aktu&#xFFFD; (*aktu&#xFFFD; (*aktu&#xFFFD; (*aktu&#xFFFD; (*aktu&#xFFFD; (*aktu&#xFFFD; (*aktu&#xFFFD; (*aktu&#xFFFD; (*aktu&#xFFFD; (*aktu&#xFFFD; (*aktu&#xFFFD; (*aktu&#xFFFD; (*aktu&#xFFFD; (*aktu&#xFFFD; (*aktu&#xFFFD; (*aktu&#xFFFD; (*aktu&#xFFFD; (*aktu&#xFFFD; (*aktu&#xFFFD; (*aktu&#xFFFD; (*aktu&#xFFFD; (*aktu&#xFFFD; (*aktu&#xFFFD; (*aktu&#xFFFD; (*aktu&#xFFFD; (*aktu&#xFFFD; (*aktu&#xFFFD; (*aktu&#xFFFD; (*aktu&#xFFFD; (*aktu&#xFFFD; (*aktu&#xFFFD; (*aktu&#xFFFD; (*aktu&#xFFFD; (*aktu&#xFFFD; (*aktu&#xFFFD; (*aktu&#xFFFD; (*aktu&#xFFFD; (*aktu&#xFFFD; (*aktu&#xFFFD; (*aktu&#xFFFD; (*aktu&#xFFFD; (*aktu&#xFFFD; (*aktu&#xFFFD; (*aktu&#xFFFD; (*aktu&#xFFFD; (*aktu&#xFFFD; (*aktu&#xFFFD; (*aktu&#xFFFD; (*aktu&#xFFFD; (*aktu&#xFFFD; (*aktu&#xFFFD; (*aktu&#xFFFD; (*aktu&#xFFFD; (*aktu&#xFFFD; (*aktu&#xFFFD; (*aktu&#xFFFD; (*aktu&#xFFFD; (*aktu&#xFFFD; (*aktu&#xFFFD; (*aktu&#xFFFD; (*aktu&#xFFFD; (*aktu&#xFFFD; (*aktu&#xFFFD; (*aktu&#xFFFD; (*aktu&#xFFFD; (*aktu&#xFFFD; (*aktu&#xFFFD; (*aktu&#xFFFD; (*aktu&#xFFFD; (*aktu&#xFFFD; (*aktu&#xFFFD; (*aktu&#xFFFD; (*aktu&#xFFFD; (*aktu&#xFFFD; (*aktu&#xFFFD; (*aktu&#xFFFD; (*aktu&#xFFFD; (*aktu&#xFFFD; (*aktu&#xFFFD; (*aktu&#xFFFD; (*aktu&#xFFFD; (*aktu&#xFFFD; (*aktu&#xFFFD; (*aktu&#xFFFD; (*aktu&#xFFFD; (*aktu&#xFFFD; (*aktu&#xFFFD; (*aktu&#xFFFD; (*aktu&#xFFFD; (*aktu&#xFFFD; (*aktu&#xFFFD; (*aktu&#xFFFD; (*aktu&#xFFFD; (*aktu&#xFFFD; (*aktu&#xFFFD; (*aktu&#xFFFD; (*aktu&#xFFFD; (*aktu&#xFFFD; (*aktu&#xFFFD; (*aktu&#xFFFD; (*aktu&#xFFFD; (*aktu&#xFFFD; (*aktu&#xFFFD; (*aktu&#xFFFD; (*aktu&#xFFFD; (*aktu&#xFFFD; (*aktu&#xFFFD; (*aktu&#xFFFD; (*aktu&#xFFFD; (*aktu&#xFFFD; (*aktu&#xFFFD; (*aktu&#xFFFD; (*aktu&#xFFFD; (*aktu&#xFFFD; (*aktu&#xFFFD; (*aktu&#xFFFD; (*aktu&#xFFFD; (*aktu&#xFFFD; (*aktu&#xFFFD; (*aktu&#xFFFD; (*aktu&#xFFFD; (*aktu&#xFFFD; (*aktu&#xFFFD; (*aktu&#xFFFD; (*aktu&#xFFFD; (*aktu&#xFFFD; (*aktu&#xFFFD; (*aktu&#xFFFD; (*aktu&#xFFFD; (*aktu&#xFFFD; (*aktu&#xFFFD; (*aktu&#xFFFD; (*aktu&#xFFFD; (*aktu&#xFFFD; (*aktu&#xFFFD; (*aktu&#xFFFD; (*aktu&#xFFFD; (*aktu&#xFFFD; (*aktu&#xFFFD; (*aktu&#xFFFD; (*aktu&#xFFFD; (*aktu&#xFFFD; (*aktu&#xFFFD; (*aktu&#xFFFD; (*aktu&#xFFFD; (*aktu&#xFFFD; (*aktu&#xFFFD; (*aktu&#xFFFD; (*aktu&#xFFFD; (*aktu&#xFFFD; (*aktu&#xFFFD; (*aktu&#xFFFD; (*aktu&#xFFFD; (*aktu&#xFFFD; (*aktu&#xFFFD; (*aktu&#xFFFD; (*aktu&#xFFFD; (*aktu&#xFFFD; (*aktu&#xFFFD; (*aktu&#xFFFD; (*aktu&#xFFFD; (*aktu&#xFFFD; (*aktu&#xFFFD; (*aktu&#xFFFD; (*aktu&#xFFFD; (*aktu&#xFFFD; (*aktu&#xFFFD; (*aktu&#xFFFD; (*aktu&#xFFFD; (*aktu&#xFFFD; (*aktu&#xFFFD; (*aktu&#xFFFD; (*aktu&#xFFFD; (*aktu&#xFFFD; (*aktu&#xFFFD; (*aktu&#xFFFD; (*aktu&#xFFFD; (*aktu&#xFFFD; (*aktu&#xFFFD; (*aktu&#xFFFD; (*aktu&#xFFFD; (*aktu&#xFFFD; (*aktu&#xFFFD; (*aktu&#xFFFD; (*aktu&#xFFFD; (*aktu&#xFFFD; (*aktu&#xFFFD; (*aktu&#xFFFD; (*aktu&#xFFFD; (*aktu&#xFFFD; (*aktu&#xFFFD; (*aktu&#xFFFD; (*aktu&#xFFFD; (*aktu&#xFFFD; (*aktu&#xFFFD; (*aktu&#xFFFD; (*aktu&#xFFFD; (*aktu&#xFFFD; (*aktu&#xFFFD; (*aktu&#xFFFD; (*aktu&#xFFFD; (*aktu&#xFFFD; (*aktu&#xFFFD; (*aktu&#xFFFD; (*aktu&#xFFFD; (*aktu&#xFFFD; (*aktu&#xFFFD; (*aktu&#xFFFD; (*aktu&#xFFFD; (*aktu&#xFFFD; (*aktu&#xFFFD; (*aktu&#xFFFD; (*aktu&#xFFFD; (*aktu&#xFFFD; (*aktu&#xFFFD; (*aktu&#xFFFD; (*aktu&#xFFFD; (*aktu&#xFFFD; (*aktu&#xFFFD; (*aktu&#xFFFD; (*aktu&#xFFFD; (*aktu&#xFFFD; (*aktu&#xFFFD; (*aktu&#xFFFD; (*aktu&#xFFFD; (*aktu&#xFFFD; (*aktu&#xFFFD; (*aktu&#xFFFD; (*aktu&#xFFFD; (*aktu&#xFFFD; (*aktu&#xFFFD; (*aktu&#xFFFD; (*aktu&#xFFFD; (*aktu&#xFFFD; (*aktu&#xFFFD; (*aktu&#xFFFD; (*aktu&#xFFFD; (*aktu&#xFFFD; (*aktu&#xFFFD; (*aktu&#xFFFD; (*aktu&#xFFFD; (*aktu&#xFFFD; (*aktu&#xFFFD; (*aktu&#xFFFD; (*aktu&#xFFFD; (*aktu&#xFFFD; (*aktu&#xFFFD; (*aktu&#xFFFD; (*aktu&#xFFFD; (*aktu&#xFFFD; (*aktu&#xFFFD; (*aktu&#xFFFD; (*aktu&#xFFFD; (*aktu&#xFFFD; (*aktu&#xFFFD; (*aktu&#xFFFD; (*aktu&#xFFFD; (*aktu&#xFFFD; (*aktu&#xFFFD; (*aktu&#xFFFD; (*aktu&#xFFFD; (*aktu&#xFFFD; (*aktu&#xFFFD; (*aktu&#xFFFD; (*aktu&#xFFFD; (*aktu&#xFFFD; (*aktu&#xFFFD; (*aktu&#xFFFD; (*aktu&#xFFFD; (*aktu&#xFFFD; (*aktu&#xFFFD; (*aktu&#xFFFD; (*aktu&#xFFFD; (*aktu&#xFFFD; (*aktu&#xFFFD; (*aktu&#xFFFD; (*aktu&#xFFFD; (*aktu&#xFFFD; (*aktu&#xFFFD; (*aktu&#xFFFD; (*aktu&#xFFFD; (*aktu&#xFFFD; (*aktu&#xFFFD; (*aktu&#xFFFD; (*aktu&#xFFFD; (*aktu&#xFFFD; (*aktu&#xFFFD; (*aktu&#xFFFD; (*aktu&#xFFFD; (*aktu&#xFFFD; (*aktu&#xFFFD; (*aktu&#xFFFD; (*aktu&#xFFFD; (*aktu&#xFFFD; (*aktu&#xFFFD; (*aktu&#xFFFD; (*aktu&#xFFFD; (*aktu&#xFFFD; (*aktu&#xFFFD; (*aktu&#xFFFD; (*aktu&#xFFFD; (*aktu&#xFFFD; (*aktu&#xFFFD; (*aktu&#xFFFD; (*aktu&#xFFFD; (*aktu&#xFFFD; (*aktu&#xFFFD; (*aktu&#xFFFD; (*aktu&#xFFFD; (*aktu&#xFFFD; (*aktu&#xFFFD; (*aktu&#xFFFD; (*aktu&#xFFFD; (*aktu&#xFFFD; (*aktu&#xFFFD; (*aktu&#xFFFD; (*aktu&#xFFFD; (*aktu&#xFFFD; (*aktu&#xFFFD; (*aktu&#xFFFD; (*aktu&#xFFFD; (*aktu&#xFFFD; (*aktu&#xFFFD; (*aktu&#xFFFD; (*aktu&#xFFFD; (*aktu&#xFFFD; (*aktu&#xFFFD; (*aktu&#xFFFD; (*aktu&#xFFFD; (*aktu&#xFFFD; (*aktu&#xFFFD; (*aktu&#xFFFD; (*aktu&#xFFFD; (*aktu&#xFFFD; (*aktu&#xFFFD; (*aktu&#xFFFD; (*aktu&#xFFFD; (*aktu&#xFFFD; (*aktu&#xFFFD; (*aktu&#xFFFD; (*aktu&#xFFFD; (*aktu&#xFFFD; (*aktu&#xFFFD; (*aktu&#xFFFD; (*aktu&#xFFFD; (*aktu&#xFFFD; (*aktu&#xFFFD; (*aktu&#xFFFD; (*aktu&#xFFFD; (*aktu&#xFFFD; (*aktu&#xFFFD; (*aktu&#xFFFD; (*aktu&#xFFFD; (*aktu&#xFFFD; (*aktu&#xFFFD; (*aktu&#xFFFD; (*aktu&#xFFFD; (*aktu&#xFFFD; (*aktu&#xFFFD; (*aktu&#xFFFD; (*aktu&#xFFFD; (*aktu&#xFFFD; (*aktu&#xFFFD; (*aktu&#xFFFD; (*aktu&#xFFFD; (*aktu&#xFFFD; (*aktu&#xFFFD; (*aktu&#xFFFD; (*aktu&#xFFFD; (*aktu&#xFFFD; (*aktu&#xFFFD; (*aktu&#xFFFD; (*aktu&#xFFFD; (*aktu&#xFFFD; (*aktu&#xFFFD; (*aktu&#xFFFD; (*aktu&#xFFFD; (*aktu&#xFFFD; (*aktu&#xFFFD; (*aktu&#xFFFD; (*aktu&#xFFFD; (*aktu&#xFFFD; (*aktu&#xFFFD; (*aktu&#xFFFD; (*aktu&#xFFFD; (*aktu&#xFFFD; (*aktu&#xFFFD; (*aktu&#xFFFD; (*aktu&#xFFFD; (*aktu&#xFFFD; (*aktu&#xFFFD; (*aktu&#xFFFD; (*aktu&#xFFFD; (*aktu&#xFFFD; (*aktu&#xFFFD; (*aktu&#xFFFD; (*aktu&#xFFFD; (*aktu&#xFFFD; (*aktu&#xFFFD; (*aktu&#xFFFD; (*aktu&#xFFFD; (*aktu&#xFFFD; (*aktu&#xFFFD; (*aktu&#xFFFD; (*aktu&#xFFFD; (*aktu&#xFFFD; (*aktu&#xFFFD; (*aktu&#xFFFD; (*aktu&#xFFFD; (*aktu&#xFFFD; (*aktu&#xFFFD; (*aktu&#xFFFD; (*aktu&#xFFFD; (*aktu&#xFFFD; (*aktu&#xFFFD; (*aktu&#xFFFD; (*aktu&#xFFFD; (*aktu&#xFFFD; (*aktu&#xFFFD; (*aktu&#xFFFD; (*aktu&#xFFFD; (*aktu&#xFFFD; (*aktu&#xFFFD; (*aktu&#xFFFD; (*aktu&#xFFFD; (*aktu&#xFFFD; (*aktu&#xFFFD; (*aktu&#xFFFD; (*aktu&#xFFFD; (*aktu&#xFFFD; (*aktu&#xFFFD; (*aktu&#xFFFD; (*aktu&#xFFFD; (*aktu&#xFFFD; (*aktu&#xFFFD; (*aktu&#xFFFD; (*aktu&#xFFFD; (*aktu&#xFFFD; (*aktu&#xFFFD; (*aktu&#xFFFD; (*aktu&#xFFFD; (*aktu&#xFFFD; (*aktu&#xFFFD; (*aktu&#xFFFD; (*aktu&#xFFFD; (*aktu&#xFFFD; (*aktu&#xFFFD; (*aktu&#xFFFD; (*aktu&#xFFFD; (*aktu&#xFFFD; (*aktu&#xFFFD; (*aktu&#xFFFD; (*aktu&#xFFFD; (*aktu&#xFFFD; (*aktu&#xFFFD; (*aktu&#xFFFD; (*aktu&#xFFFD; (*aktu&#xFFFD; (*aktu&#xFFFD; (*aktu&#xFFFD; (*aktu&#xFFFD; (*aktu&#xFFFD; (*aktu&#xFFFD; (*aktu&#xFFFD; (*aktu&#xFFFD; (*aktu&#xFFFD; (*aktu&#xFFFD; (*aktu&#xFFFD; (*aktu&#xFFFD; (*aktu&#xFFFD; (*aktu&#xFFFD; (*aktu&#xFFFD; (*aktu&#xFFFD; (*aktu&#xFFFD; (*aktu&#xFFFD; (*aktu&#xFFFD; (*aktu&#xFFFD; (*aktu&#xFFFD; (*aktu&#xFFFD; (*aktu&#xFFFD; (*aktu&#xFFFD; (*aktu&#xFFFD; (*aktu&#xFFFD; (*aktu&#xFFFD; (*aktu&#xFFFD; (*aktu&#xFFFD; (*aktu&#xFFFD; (*aktu&#xFFFD; (*aktu&#xFFFD; (*aktu&#xFFFD; (*aktu&#xFFFD; (*aktu&#xFFFD; (*aktu&#xFFFD; (*aktu&#xFFFD; (*aktu&#xFFFD; (*aktu&#xFFFD; (*aktu&#xFFFD; (*aktu&#xFFFD; (*aktu&#xFFFD; (*aktu&#xFFFD; (*aktu&#xFFFD; (*aktu&#xFFFD; (*aktu&#xFFFD; (*aktu&#xFFFD; (*aktu&#xFFFD; (*aktu&#xFFFD; (*aktu&#xFFFD; (*aktu&#xFFFD; (*aktu&#xFFFD; (*aktu&#xFFFD; (*aktu&#xFFFD; (*aktu&#xFFFD; (*aktu&#xFFFD; (*aktu&#xFFFD; (*aktu&#xFFFD; (*aktu&#xFFFD; (*aktu&#xFFFD; (*aktu&#xFFFD; (*aktu&#xFFFD; (*aktu&#xFFFD; (*aktu&#xFFFD; (*aktu&#xFFFD; (*aktu&#xFFFD; (*aktu&#xFFFD; (*aktu&#xFFFD; (*aktu&#xFFFD; (*aktu&#xFFFD; (*aktu&#xFFFD; (*aktu&#xFFFD; (*aktu&#xFFFD; (*aktu&#xFFFD; (*aktu&#xFFFD; (*aktu&#xFFFD; (*aktu&#xFFFD; (*aktu&#xFFFD; (*aktu&#xFFFD; (*aktu&#xFFFD; (*aktu&#xFFFD; (*aktu&#xFFFD; (*aktu&#xFFFD; (*aktu&#xFFFD; (*aktu&#xFFFD; (*aktu&#xFFFD; (*aktu&#xFFFD; (*aktu&#xFFFD; (*aktu&#xFFFD; (*aktu&#xFFFD; (*aktu&#xFFFD; (*aktu&#xFFFD; (*aktu&#xFFFD; (*aktu&#xFFFD; (*aktu&#xFFFD; (*aktu&#xFFFD; (*aktu&#xFFFD; (*aktu&#xFFFD; (*aktu&#xFFFD; (*aktu&#xFFFD; (*aktu&#xFFFD; (*aktu&#xFFFD; (*aktu&#xFFFD; (*aktu&#xFFFD; (*aktu&#xFFFD; (*aktu&#xFFFD; (*aktu&#xFFFD; (*aktu&#xFFFD; (*aktu&#xFFFD; (*aktu&#xFFFD; (*aktu&#xFFFD; (*aktu&#xFFFD; (*aktu&#xFFFD; (*aktu&#xFFFD; (*aktu&#xFFFD; (*aktu&#xFFFD; (*aktu&#xFFFD; (*aktu&#xFFFD; (*aktu&#xFFFD; (*aktu&#xFFFD; (*aktu&#xFFFD; (*aktu&#xFFFD; (*aktu&#xFFFD; (*aktu&#xFFFD; (*aktu&#xFFFD; (*aktu&#xFFFD; (*aktu&#xFFFD; (*aktu&#xFFFD; (*aktu&#xFFFD; (*aktu&#xFFFD; (*aktu&#xFFFD; (*aktu&#xFFFD; (*aktu&#xFFFD; (*aktu&#xFFFD; (*aktu&#xFFFD; (*aktu&#xFFFD; (*aktu&#xFFFD; (*aktu&#xFFFD; (*aktu&#xFFFD; (*aktu&#xFFFD; (*aktu&#xFFFD; (*aktu&#xFFFD; (*aktu&#xFFFD; (*aktu&#xFFFD; (*aktu&#xFFFD; (*aktu&#xFFFD; (*aktu&#xFFFD; (*aktu&#xFFFD; (*aktu&#xFFFD; (*aktu&#xFFFD; (*aktu&#xFFFD; (*aktu&#xFFFD; (*aktu&#xFFFD; (*aktu&#xFFFD; (*aktu&#xFFFD; (*aktu&#xFFFD; (*aktu&#xFFFD; (*aktu&#xFFFD; (*aktu&#xFFFD; (*aktu&#xFFFD; (*aktu&#xFFFD; (*aktu&#xFFFD; (*aktu&#xFFFD; (*aktu&#xFFFD; (*aktu&#xFFFD; (*aktu&#xFFFD; (*aktu&#xFFFD; (*aktu&#xFFFD; (*aktu&#xFFFD; (*aktu&#xFFFD; (*aktu&#xFFFD; (*aktu&#xFFFD; (*aktu&#xFFFD; (*aktu&#xFFFD; (*aktu&#xFFFD; (*aktu&#xFFFD; (*aktu&#xFFFD; (*aktu&#xFFFD; (*aktu&#xFFFD; (*aktu&#xFFFD; (*aktu&#xFFFD; (*aktu&#xFFFD; (*aktu&#xFFFD; (*aktu&#xFFFD; (*aktu&#xFFFD; (*aktu&#xFFFD; (*aktu&#xFFFD; (*aktu&#xFFFD; (*aktu&#xFFFD; (*aktu&#xFFFD; (*aktu&#xFFFD; (*aktu&#xFFFD; (*aktu&#xFFFD; (*aktu&#xFFFD; (*aktu&#xFFFD; (*aktu&#xFFFD; (*aktu&#xFFFD; (*aktu&#xFFFD; (*aktu&#xFFFD; (*aktu&#xFFFD; (*aktu&#xFFFD; (*aktu&#xFFFD; (*aktu&#xFFFD; (*aktu&#xFFFD; (*aktu&#xFFFD; (*aktu&#xFFFD; (*aktu&#xFFFD; (*aktu&#xFFFD; (*aktu&#xFFFD; (*aktu&#xFFFD; (*aktu&#xFFFD; (*aktu&#xFFFD; (*aktu&#xFFFD; (*aktu&#xFFFD; (*aktu&#xFFFD; (*aktu&#xFFFD; (*aktu&#xFFFD; (*aktu&#xFFFD; (*aktu&#xFFFD; (*aktu&#xFFFD; (*aktu&#xFFFD; (*aktu&#xFFFD; (*aktu&#xFFFD; (*aktu&#xFFFD; (*aktu&#xFFFD; (*aktu&#xFFFD; (*aktu&#xFFFD; (*aktu&#xFFFD; (*aktu&#xFFFD; (*aktu&#xFFFD; (*aktu&#xFFFD; (*aktu&#xFFFD; (*aktu&#xFFFD; (*aktu&#xFFFD; (*aktu&#xFFFD; (*aktu&#xFFFD; (*aktu&#xFFFD; (*aktu&#xFFFD; (*aktu&#xFFFD; (*aktu&#xFFFD; (*aktu&#xFFFD; (*aktu&#xFFFD; (*aktu&#xFFFD; (*aktu&#xFFFD; (*aktu&#xFFFD; (*aktu&#xFFFD; (*aktu&#xFFFD; (*aktu&#xFFFD; (*aktu&#xFFFD; (*aktu&#xFFFD; (*aktu&#xFFFD; (*aktu&#xFFFD; (*aktu&#xFFFD; (*aktu&#xFFFD; (*aktu&#xFFFD; (*aktu&#xFFFD; (*aktu&#xFFFD; (*aktu&#xFFFD; (*aktu&#xFFFD; (*aktu&#xFFFD; (*aktu&#xFFFD; (*aktu&#xFFFD; (*aktu&#xFFFD; (*aktu&#xFFFD; (*aktu&#xFFFD; (*aktu&#xFFFD; (*aktu&#xFFFD; (*aktu&#xFFFD; (*aktu&#xFFFD; (*aktu&#xFFFD; (*aktu&#xFFFD; (*aktu&#xFFFD; (*aktu&#xFFFD; (*aktu&#xFFFD; (*aktu&#xFFFD; (*aktu&#xFFFD; (*aktu&#xFFFD; (*aktu&#xFFFD; (*aktu&#xFFFD; (*aktu&#xFFFD; (*aktu&#xFFFD; (*aktu&#xFFFD; (*aktu&#xFFFD; (*aktu&#xFFFD; (*aktu&#xFFFD; (*aktu&#xFFFD; (*aktu&#xFFFD; (*aktu&#xFFFD; (*aktu&#xFFFD; (*aktu&#xFFFD; (*aktu&#xFFFD; (*aktu&#xFFFD; (*aktu&#xFFFD; (*aktu&#xFFFD; (*aktu&#xFFFD; (*aktu&#xFFFD; (*aktu&#xFFFD; (*aktu&#xFFFD; (*aktu&#xFFFD; (*aktu&#xFFFD; (*aktu&#xFFFD; (*aktu&#xFFFD; (*aktu&#xFFFD; (*aktu&#xFFFD; (*aktu&#xFFFD; (*aktu&#xFFFD; (*aktu&#xFFFD; (*aktu&#xFFFD; (*aktu&#xFFFD; (*aktu&#xFFFD; (*aktu&#xFFFD; (*aktu&#xFFFD; (*aktu&#xFFFD; (*aktu&#xFFFD; (*aktu&#xFFFD; (*aktu&#xFFFD; (*aktu&#xFFFD; (*aktu&#xFFFD; (*aktu&#xFFFD; (*aktu&#xFFFD; (*aktu&#xFFFD; (*aktu&#xFFFD; (*aktu&#xFFFD; (*aktu&#xFFFD; (*aktu&#xFFFD; (*aktu&#xFFFD; (*aktu&#xFFFD; (*aktu&#xFFFD; (*aktu&#xFFFD; (*aktu&#xFFFD; (*aktu&#xFFFD; (*aktu&#xFFFD; (*aktu&#xFFFD; (*aktu&#xFFFD; (*aktu&#xFFFD; (*aktu&#xFFFD; (*aktu&#xFFFD; (*aktu&#xFFFD; (*aktu&#xFFFD; (*aktu&#xFFFD; (*aktu&#xFFFD; (*aktu&#xFFFD; (*aktu&#xFFFD; (*aktu&#xFFFD; (*aktu&#xFFFD; (*aktu&#xFFFD; (*aktu&#xFFFD; (*aktu&#xFFFD; (*aktu&#xFFFD; (*aktu&#xFFFD; (*aktu&#xFFFD; (*aktu&#xFFFD; (*aktu&#xFFFD; (*aktu&#xFFFD; (*aktu&#xFFFD; (*aktu&#xFFFD; (*aktu&#xFFFD; (*aktu&#xFFFD; (*aktu&#xFFFD; (*aktu&#xFFFD; (*aktu&#xFFFD; (*aktu&#xFFFD; (*aktu&#xFFFD; (*aktu&#xFFFD; (*aktu&#xFFFD; (*aktu&#xFFFD; (*aktu&#xFFFD; (*aktu&#xFFFD; (*aktu&#xFFFD; (*aktu&#xFFFD; (*aktu&#xFFFD; (*aktu&#xFFFD; (*aktu&#xFFFD; (*aktu&#xFFFD; (*aktu&#xFFFD; (*aktu&#xFFFD; (*aktu&#xFFFD; (*aktu&#xFFFD; (*aktu&#xFFFD; (*aktu&#xFFFD; (*aktu&#xFFFD; (*aktu&#xFFFD; (*aktu&#xFFFD; (*aktu&#xFFFD; (*aktu&#xFFFD; (*aktu&#xFFFD; (*aktu&#xFFFD; (*aktu&#xFFFD; (*aktu&#xFFFD; (*aktu&#xFFFD; (*aktu&#xFFFD; (*aktu&#xFFFD; (*aktu&#xFFFD; (*aktu&#xFFFD; (*aktu&#xFFFD; (*aktu&#xFFFD; (*aktu&#xFFFD; (*aktu&#xFFFD; (*aktu&#xFFFD; (*aktu&#xFFFD; (*aktu&#xFFFD; (*aktu&#xFFFD; (*aktu&#xFFFD; (*aktu&#xFFFD; (*aktu&#xFFFD; (*aktu&#xFFFD; (*aktu&#xFFFD; (*aktu&#xFFFD; (*aktu&#xFFFD; (*aktu&#xFFFD; (*aktu&#xFFFD; (*aktu&#xFFFD; (*aktu&#xFFFD; (*aktu&#xFFFD; (*aktu&#xFFFD; (*aktu&#xFFFD; (*aktu&#xFFFD; (*aktu&#xFFFD; (*aktu&#xFFFD; (*aktu&#xFFFD; (*aktu&#xFFFD; (*aktu&#xFFFD; (*aktu&#xFFFD; (*aktu&#xFFFD; (*aktu&#xFFFD; (*aktu&#xFFFD; (*aktu&#xFFFD; (*aktu&#xFFFD; (*aktu&#xFFFD; (*aktu&#xFFFD; (*aktu&#xFFFD; (*aktu&#xFFFD; (*aktu&#xFFFD; (*aktu&#xFFFD; (*aktu&#xFFFD; (*aktu&#xFFFD; (*aktu&#xFFFD; (*aktu&#xFFFD; (*aktu&#xFFFD; (*aktu&#xFFFD; (*aktu&#xFFFD; (*aktu&#xFFFD; (*aktu&#xFFFD; (*aktu&#xFFFD; (*aktu&#xFFFD; (*aktu&#xFFFD; (*aktu&#xFFFD; (*aktu&#xFFFD; (*aktu&#xFFFD; (*aktu&#xFFFD; (*aktu&#xFFFD; (*aktu&#xFFFD; (*aktu&#xFFFD; (*aktu&#xFFFD; (*aktu&#xFFFD; (*aktu&#xFFFD; (*aktu&#xFFFD; (*aktu&#xFFFD; (*aktu&#xFFFD; (*aktu&#xFFFD; (*aktu&#xFFFD; (*aktu&#xFFFD; (*aktu&#xFFFD; (*aktu&#xFFFD; (*aktu&#xFFFD; (*aktu&#xFFFD; (*aktu&#xFFFD; (*aktu&#xFFFD; (*aktu&#xFFFD; (*aktu&#xFFFD; (*aktu&#xFFFD; (*aktu&#xFFFD; (*aktu&#xFFFD; (*aktu&#xFFFD; (*aktu&#xFFFD; (*aktu&#xFFFD; (*aktu&#xFFFD; (*aktu&#xFFFD; (*aktu&#xFFFD; (*aktu&#xFFFD; (*aktu&#xFFFD; (*aktu&#xFFFD; (*aktu&#xFFFD; (*aktu&#xFFFD; (*aktu&#xFFFD; (*aktu&#xFFFD; (*aktu&#xFFFD; (*aktu&#xFFFD; (*aktu&#xFFFD; (*aktu&#xFFFD; (*aktu&#xFFFD; (*aktu&#xFFFD; (*aktu&#xFFFD; (*aktu&#xFFFD; (*aktu&#xFFFD; (*aktu&#xFFFD; (*aktu&#xFFFD; (*aktu&#xFFFD; (*aktu&#xFFFD; (*aktu&#xFFFD; (*aktu&#xFFFD; (*aktu&#xFFFD; (*aktu&#xFFFD; (*aktu&#xFFFD; (*aktu&#xFFFD; (*aktu&#xFFFD; (*aktu&#xFFFD; (*aktu&#xFFFD; (*aktu&#xFFFD; (*aktu&#xFFFD; (*aktu&#xFFFD; (*aktu&#xFFFD; (*aktu&#xFFFD; (*aktu&#xFFFD; (*aktu&#xFFFD; (*aktu&#xFFFD; (*aktu&#xFFFD; (*aktu&#xFFFD; (*aktu&#xFFFD; (*aktu&#xFFFD; (*aktu&#xFFFD; (*aktu&#xFFFD; (*aktu&#xFFFD; (*aktu&#xFFFD; (*aktu&#xFFFD; (*aktu&#xFFFD; (*aktu&#xFFFD; (*aktu&#xFFFD; (*aktu&#xFFFD; (*aktu&#xFFFD; (*aktu&#xFFFD; (*aktu&#xFFFD; (*aktu&#xFFFD; (*aktu&#xFFFD; (*aktu&#xFFFD; (*aktu&#xFFFD; (*aktu&#xFFFD; (*aktu&#xFFFD; (*aktu&#xFFFD; (*aktu&#xFFFD; (*aktu&#xFFFD; (*aktu&#xFFFD; (*aktu&#xFFFD; (*aktu&#xFFFD; (*aktu&#xFFFD; (*aktu&#xFFFD; (*aktu&#xFFFD; (*aktu&#xFFFD; (*aktu&#xFFFD; (*aktu&#xFFFD; (*aktu&#xFFFD; (*aktu&#xFFFD; (*aktu&#xFFFD; (*aktu&#xFFFD; (*aktu&#xFFFD; (*aktu&#xFFFD; (*aktu&#xFFFD; (*aktu&#xFFFD; (*aktu&#xFFFD; (*aktu&#xFFFD; (*aktu&#xFFFD; (*aktu&#xFFFD; (*aktu&#xFFFD; (*aktu&#xFFFD; (*aktu&#xFFFD; (*aktu&#xFFFD; (*aktu&#xFFFD; (*aktu&#xFFFD; (*aktu&#xFFFD; (*aktu&#xFFFD; (*aktu&#xFFFD; (*aktu&#xFFFD; (*aktu&#xFFFD; (*aktu&#xFFFD; (*aktu&#xFFFD; (*aktu&#xFFFD; (*aktu&#xFFFD; (*aktu&#xFFFD; (*aktu&#xFFFD; (*aktu&#xFFFD; (*aktu&#xFFFD; (*aktu&#xFFFD; (*aktu&#xFFFD; (*aktu&#xFFFD; (*aktu&#xFFFD; (*aktu&#xFFFD; (*aktu&#xFFFD; (*aktu&#xFFFD; (*aktu&#xFFFD; (*aktu&#xFFFD; (*aktu&#xFFFD; (*aktu&#xFFFD; (*aktu&#xFFFD; (*aktu&#xFFFD; (*aktu&#xFFFD; (*aktu&#xFFFD; (*aktu&#xFFFD; (*aktu&#xFFFD; (*aktu&#xFFFD; (*aktu&#xFFFD; (*aktu&#xFFFD; (*aktu&#xFFFD; (*aktu&#xFFFD; (*aktu&#xFFFD; (*aktu&#xFFFD; (*aktu&#xFFFD; (*aktu&#xFFFD; (*aktu&#xFFFD; (*aktu&#xFFFD; (*aktu&#xFFFD; (*aktu&#xFFFD; (*aktu&#xFFFD; (*aktu&#xFFFD; (*aktu&#xFFFD; (*aktu&#xFFFD; (*aktu&#xFFFD; (*aktu&#xFFFD; (*aktu&#xFFFD; (*aktu&#xFFFD; (*aktu&#xFFFD; (*aktu&#xFFFD; (*aktu&#xFFFD; (*aktu&#xFFFD; (*aktu&#xFFFD; (*aktu&#xFFFD; (*aktu&#xFFFD; (*aktu&#xFFFD; (*aktu&#xFFFD; (*aktu&#xFFFD; (*aktu&#xFFFD; (*aktu&#xFFFD; (*aktu&#xFFFD; (*aktu&#xFFFD; (*aktu&#xFFFD; (*aktu&#xFFFD; (*aktu&#xFFFD; (*aktu&#xFFFD; (*aktu&#xFFFD; (*aktu&#xFFFD; (*aktu&#xFFFD; (*aktu&#xFFFD; (*aktu&#xFFFD; (*aktu&#xFFFD; (*aktu&#xFFFD; (*aktu&#xFFFD; (*aktu&#xFFFD; (*aktu&#xFFFD; (*aktu&#xFFFD; (*aktu&#xFFFD; (*aktu&#xFFFD; (*aktu&#xFFFD; (*aktu&#xFFFD; (*aktu&#xFFFD; (*aktu&#xFFFD; (*aktu&#xFFFD; (*aktu&#xFFFD; (*aktu&#xFFFD; (*aktu&#xFFFD; (*aktu&#xFFFD; (*aktu&#xFFFD; (*aktu&#xFFFD; (*aktu&#xFFFD; (*aktu&#xFFFD; (*aktu&#xFFFD; (*aktu&#xFFFD; (*aktu&#xFFFD; (*aktu&#xFFFD; (*aktu&#xFFFD; (*aktu&#xFFFD; (*aktu&#xFFFD; (*aktu&#xFFFD; (*aktu&#xFFFD; (*aktu&#xFFFD; (*aktu&#xFFFD; (*aktu&#xFFFD; (*aktu&#xFFFD; (*aktu&#xFFFD; (*aktu&#xFFFD; (*aktu&#xFFFD; (*aktu&#xFFFD; (*aktu&#xFFFD; (*aktu&#xFFFD; (*aktu&#xFFFD; (*aktu&#xFFFD; (*aktu&#xFFFD; (*aktu&#xFFFD; (*aktu&#xFFFD; (*aktu&#xFFFD; (*aktu&#xFFFD; (*aktu&#xFFFD; (*aktu&#xFFFD; (*aktu&#xFFFD; (*aktu&#xFFFD; (*aktu&#xFFFD; (*aktu&#xFFFD; (*aktu&#xFFFD; (*aktu&#xFFFD; (*aktu&#xFFFD; (*aktu&#xFFFD; (*aktu&#xFFFD; (*aktu&#xFFFD; (*aktu&#xFFFD; (*aktu&#xFFFD; (*aktu&#xFFFD; (*aktu&#xFFFD; (*aktu&#xFFFD; (*aktu&#xFFFD; (*aktu&#xFFFD; (*aktu&#xFFFD; (*aktu&#xFFFD; (*aktu&#xFFFD; (*aktu&#xFFFD; (*aktu&#xFFFD; (*aktu&#xFFFD; (*aktu&#xFFFD; (*aktu&#xFFFD; (*aktu&#xFFFD; (*aktu&#xFFFD; (*aktu&#xFFFD; (*aktu&#xFFFD; (*aktu&#xFFFD; (*aktu&#xFFFD; (*aktu&#xFFFD; (*aktu&#xFFFD; (*aktu&#xFFFD; (*aktu&#xFFFD; (*aktu&#xFFFD; (*aktu&#xFFFD; (*aktu&#xFFFD; (*aktu&#xFFFD; (*aktu&#xFFFD; (*aktu&#xFFFD; (*aktu&#xFFFD; (*aktu&#xFFFD; (*aktu&#xFFFD; (*aktu&#xFFFD; (*aktu&#xFFFD; (*aktu&#xFFFD; (*aktu&#xFFFD; (*aktu&#xFFFD; (*aktu&#xFFFD; (*aktu&#xFFFD; (*aktu&#xFFFD; (*aktu&#xFFFD; (*aktu&#xFFFD; (*aktu&#xFFFD; (*aktu&#xFFFD; (*aktu&#xFFFD; (*aktu&#xFFFD; (*aktu&#xFFFD; (*aktu&#xFFFD; (*aktu&#xFFFD; (*aktu&#xFFFD; (*aktu&#xFFFD; (*aktu&#xFFFD; (*aktu&#xFFFD; (*aktu&#xFFFD; (*aktu&#xFFFD; (*aktu&#xFFFD; (*aktu&#xFFFD; (*aktu&#xFFFD; (*aktu&#xFFFD; (*aktu&#xFFFD; (*aktu&#xFFFD; (*aktu&#xFFFD; (*aktu&#xFFFD; (*aktu&#xFFFD; (*aktu&#xFFFD; (*aktu&#xFFFD; (*aktu&#xFFFD; (*aktu&#xFFFD; (*aktu&#xFFFD; (*aktu&#xFFFD; (*aktu&#xFFFD; (*aktu&#xFFFD; (*aktu&#xFFFD; (*aktu&#xFFFD; (*aktu&#xFFFD; (*aktu&#xFFFD; (*aktu&#xFFFD; (*aktu&#xFFFD; (*aktu&#xFFFD; (*aktu&#xFFFD; (*aktu&#xFFFD; (*aktu&#xFFFD; (*aktu&#xFFFD; (*aktu&#xFFFD; (*aktu&#xFFFD; (*aktu&#xFFFD; (*aktu&#xFFFD; (*aktu&#xFFFD; (*aktu&#xFFFD; (*aktu&#xFFFD; (*aktu&#xFFFD; (*aktu&#xFFFD; (*aktu&#xFFFD; (*aktu&#xFFFD; (*aktu&#xFFFD; (*aktu&#xFFFD; (*aktu&#xFFFD; (*aktu&#xFFFD; (*aktu&#xFFFD; (*aktu&#xFFFD; (*aktu&#xFFFD; (*aktu&#xFFFD; (*aktu&#xFFFD; (*aktu&#xFFFD; (*aktu&#xFFFD; (*aktu&#xFFFD; (*aktu&#xFFFD; (*aktu&#xFFFD; (*aktu&#xFFFD; (*aktu&#xFFFD; (*aktu&#xFFFD; (*aktu&#xFFFD; (*aktu&#xFFFD; (*aktu&#xFFFD; (*aktu&#xFFFD; (*aktu&#xFFFD; (*aktu&#xFFFD; (*aktu&#xFFFD; (*aktu&#xFFFD; (*aktu&#xFFFD; (*aktu&#xFFFD; (*aktu&#xFFFD; (*aktu&#xFFFD; (*aktu&#xFFFD; (*aktu&#xFFFD; (*aktu&#xFFFD; (*aktu&#xFFFD; (*aktu&#xFFFD; (*aktu&#xFFFD; (*aktu&#xFFFD; (*aktu&#xFFFD; (*aktu&#xFFFD; (*aktu&#xFFFD; (*aktu&#xFFFD; (*aktu&#xFFFD; (*aktu&#xFFFD; (*aktu&#xFFFD; (*aktu&#xFFFD; (*aktu&#xFFFD; (*aktu&#xFFFD; (*aktu&#xFFFD; (*aktu&#xFFFD; (*aktu&#xFFFD; (*aktu&#xFFFD; (*aktu&#xFFFD; (*aktu&#xFFFD; (*aktu&#xFFFD; (*aktu&#xFFFD; (*aktu&#xFFFD; (*aktu&#xFFFD; (*aktu&#xFFFD; (*aktu&#xFFFD; (*aktu&#xFFFD; (*aktu&#xFFFD; (*aktu&#xFFFD; (*aktu&#xFFFD; (*aktu&#xFFFD; (*aktu&#xFFFD; (*aktu&#xFFFD; (*aktu&#xFFFD; (*aktu&#xFFFD; (*aktu&#xFFFD; (*aktu&#xFFFD; (*aktu&#xFFFD; (*aktu&#xFFFD; (*aktu&#xFFFD; (*aktu&#xFFFD; (*aktu&#xFFFD; (*aktu&#xFFFD; (*aktu&#xFFFD; (*aktu&#xFFFD; (*aktu&#xFFFD; (*aktu&#xFFFD; (*aktu&#xFFFD; (*aktu&#xFFFD; (*aktu&#xFFFD; (*aktu&#xFFFD; (*aktu&#xFFFD; (*aktu&#xFFFD; (*aktu&#xFFFD; (*aktu&#xFFFD; (*aktu&#xFFFD; (*aktu&#xFFFD; (*aktu&#xFFFD; (*aktu&#xFFFD; (*aktu&#xFFFD; (*aktu&#xFFFD; (*aktu&#xFFFD; (*aktu&#xFFFD; (*aktu&#xFFFD; (*aktu&#xFFFD; (*aktu&#xFFFD; (*aktu&#xFFFD; (*aktu&#xFFFD; (*aktu&#xFFFD; (*aktu&#xFFFD; (*aktu&#xFFFD; (*aktu&#xFFFD; (*aktu&#xFFFD; (*aktu&#xFFFD; (*aktu&#xFFFD; (*aktu&#xFFFD; (*aktu&#xFFFD; (*aktu&#xFFFD; (*aktu&#xFFFD; (*aktu&#xFFFD; (*aktu&#xFFFD; (*aktu&#xFFFD; (*aktu&#xFFFD; (*aktu&#xFFFD; (*aktu&#xFFFD; (*aktu&#xFFFD; (*aktu&#xFFFD; (*aktu&#xFFFD; (*aktu&#xFFFD; (*aktu&#xFFFD; (*aktu&#xFFFD; (*aktu&#xFFFD; (*aktu&#xFFFD; (*aktu&#xFFFD; (*aktu&#xFFFD; (*aktu&#xFFFD; (*aktu&#xFFFD; (*aktu&#xFFFD; (*aktu&#xFFFD; (*aktu&#xFFFD; (*aktu&#xFFFD; (*aktu&#xFFFD; (*aktu&#xFFFD; (*aktu&#xFFFD; (*aktu&#xFFFD; (*aktu&#xFFFD; (*aktu&#xFFFD; (*aktu&#xFFFD; (*aktu&#xFFFD; (*aktu&#xFFFD; (*aktu&#xFFFD; (*aktu&#xFFFD; (*aktu&#xFFFD; (*aktu&#xFFFD; (*aktu&#xFFFD; (*aktu&#xFFFD; (*aktu&#xFFFD; (*aktu&#xFFFD; (*aktu&#xFFFD; (*aktu&#xFFFD; (*aktu&#xFFFD; (*aktu&#xFFFD; (*aktu&#xFFFD; (*aktu&#xFFFD; (*aktu&#xFFFD; (*aktu&#xFFFD; (*aktu&#xFFFD; (*aktu&#xFFFD; (*aktu&#xFFFD; (*aktu&#xFFFD; (*aktu&#xFFFD; (*aktu&#xFFFD; (*aktu&#xFFFD; (*aktu&#xFFFD; (*aktu&#xFFFD; (*aktu&#xFFFD; (*aktu&#xFFFD; (*aktu&#xFFFD; (*aktu&#xFFFD; (*aktu&#xFFFD; (*aktu&#xFFFD; (*aktu&#xFFFD; (*aktu&#xFFFD; (*aktu&#xFFFD; (*aktu&#xFFFD; (*aktu&#xFFFD; (*aktu&#xFFFD; (*aktu&#xFFFD; (*aktu&#xFFFD; (*aktu&#xFFFD; (*aktu&#xFFFD; (*aktu&#xFFFD; (*aktu&#xFFFD; (*aktu&#xFFFD; (*aktu&#xFFFD; (*aktu&#xFFFD; (*aktu&#xFFFD; (*aktu&#xFFFD; (*aktu&#xFFFD; (*aktu&#xFFFD; (*aktu&#xFFFD; (*aktu&#xFFFD; (*aktu&#xFFFD; (*aktu&#xFFFD; (*aktu&#xFFFD; (*aktu&#xFFFD; (*aktu&#xFFFD; (*aktu&#xFFFD; (*aktu&#xFFFD; (*aktu&#xFFFD; (*aktu&#xFFFD; (*aktu&#xFFFD; (*aktu&#xFFFD; (*aktu&#xFFFD; (*aktu&#xFFFD; (*aktu&#xFFFD; (*aktu&#xFFFD; (*aktu&#xFFFD; (*aktu&#xFFFD; (*aktu&#xFFFD; (*aktu&#xFFFD; (*aktu&#xFFFD; (*aktu&#xFFFD; (*aktu&#xFFFD; (*aktu&#xFFFD; (*aktu&#xFFFD; (*aktu&#xFFFD; (*aktu&#xFFFD; (*aktu&#xFFFD; (*aktu&#xFFFD; (*aktu&#xFFFD; (*aktu&#xFFFD; (*aktu&#xFFFD; (*aktu&#xFFFD; (*aktu&#xFFFD; (*aktu&#xFFFD; (*aktu&#xFFFD; (*aktu&#xFFFD; (*aktu&#xFFFD; (*aktu&#xFFFD; (*aktu&#xFFFD; (*aktu&#xFFFD; (*aktu&#xFFFD; (*aktu&#xFFFD; (*aktu&#xFFFD; (*aktu&#xFFFD; (*aktu&#xFFFD; (*aktu&#xFFFD; (*aktu&#xFFFD; (*aktu&#xFFFD; (*aktu&#xFFFD; (*aktu&#xFFFD; (*aktu&#xFFFD; (*aktu&#xFFFD; (*aktu&#xFFFD; (*aktu&#xFFFD; (*aktu&#xFFFD; (*aktu&#xFFFD; (*aktu&#xFFFD; (*aktu&#xFFFD; (*aktu&#xFFFD; (*aktu&#xFFFD; (*aktu&#xFFFD; (*aktu&#xFFFD; (*aktu&#xFFFD; (*aktu&#xFFFD; (*aktu&#xFFFD; (*aktu&#xFFFD; (*aktu&#xFFFD; (*aktu&#xFFFD; (*aktu&#xFFFD; (*aktu&#xFFFD; (*aktu&#xFFFD; (*aktu&#xFFFD; (*aktu&#xFFFD; (*aktu&#xFFFD; (*aktu&#xFFFD; (*aktu&#xFFFD; (*aktu&#xFFFD; (*aktu&#xFFFD; (*aktu&#xFFFD; (*aktu&#xFFFD; (*aktu&#xFFFD; (*aktu&#xFFFD; (*aktu&#xFFFD; (*aktu&#xFFFD; (*aktu&#xFFFD; (*aktu&#xFFFD; (*aktu&#xFFFD; (*aktu&#xFFFD; (*aktu&#xFFFD; (*aktu&#xFFFD; (*aktu&#xFFFD; (*aktu&#xFFFD; (*aktu&#xFFFD; (*aktu&#xFFFD; (*aktu&#xFFFD; (*aktu&#xFFFD; (*aktu&#xFFFD; (*aktu&#xFFFD; (*aktu&#xFFFD; (*aktu&#xFFFD; (*aktu&#xFFFD; (*aktu&#xFFFD; (*aktu&#xFFFD; (*aktu&#xFFFD; (*aktu&#xFFFD; (*aktu&#xFFFD; (*aktu&#xFFFD; (*aktu&#xFFFD; (*aktu&#xFFFD; (*aktu&#xFFFD; (*aktu&#xFFFD; (*aktu&#xFFFD; (*aktu&#xFFFD; (*aktu&#xFFFD; (*aktu&#xFFFD; (*aktu&#xFFFD; (*aktu&#xFFFD; (*aktu&#xFFFD; (*aktu&#xFFFD; (*aktu&#xFFFD; (*aktu&#xFFFD; (*aktu&#xFFFD; (*aktu&#xFFFD; (*aktu&#xFFFD; (*aktu&#xFFFD; (*aktu&#xFFFD; (*aktu&#xFFFD; (*aktu&#xFFFD; (*aktu&#xFFFD; (*aktu&#xFFFD; (*aktu&#xFFFD; (*aktu&#xFFFD; (*aktu&#xFFFD; (*aktu&#xFFFD; (*aktu&#xFFFD; (*aktu&#xFFFD; (*aktu&#xFFFD; (*aktu&#xFFFD; (*aktu&#xFFFD; (*aktu&#xFFFD; (*aktu&#xFFFD; (*aktu&#xFFFD; (*aktu&#xFFFD; (*aktu&#xFFFD; (*aktu&#xFFFD; (*aktu&#xFFFD; (*aktu&#xFFFD; (*aktu&#xFFFD; (*aktu&#xFFFD; (*aktu&#xFFFD; (*aktu&#xFFFD; (*aktu&#xFFFD; (*aktu&#xFFFD; (*aktu&#xFFFD; (*aktu&#xFFFD; (*aktu&#xFFFD; (*aktu&#xFFFD; (*aktu&#xFFFD; (*aktu&#xFFFD; (*aktu&#xFFFD; (*aktu&#xFFFD; (*aktu&#xFFFD; (*aktu&#xFFFD; (*aktu&#xFFFD; (*aktu&#xFFFD; (*aktu&#xFFFD; (*aktu&#xFFFD; (*aktu&#xFFFD; (*aktu&#xFFFD; (*aktu&#xFFFD; (*aktu&#xFFFD; (*aktu&#xFFFD; (*aktu&#xFFFD; (*aktu&#xFFFD; (*aktu&#xFFFD; (*aktu&#xFFFD; (*aktu&#xFFFD; (*aktu&#xFFFD; (*aktu&#xFFFD; (*aktu&#xFFFD; (*aktu&#xFFFD; (*aktu&#xFFFD; (*aktu&#xFFFD; (*aktu&#xFFFD; (*aktu&#xFFFD; (*aktu&#xFFFD; (*aktu&#xFFFD; (*aktu&#xFFFD; (*aktu&#xFFFD; (*aktu&#xFFFD; (*aktu&#xFFFD; (*aktu&#xFFFD; (*aktu&#xFFFD; (*aktu&#xFFFD; (*aktu&#xFFFD; (*aktu&#xFFFD; (*aktu&#xFFFD; (*aktu&#xFFFD; (*aktu&#xFFFD; (*aktu&#xFFFD; (*aktu&#xFFFD; (*aktu&#xFFFD; (*aktu&#xFFFD; (*aktu&#xFFFD; (*aktu&#xFFFD; (*aktu&#xFFFD; (*aktu&#xFFFD; (*aktu&#xFFFD; (*aktu&#xFFFD; (*aktu&#xFFFD; (*aktu&#xFFFD; (*aktu&#xFFFD; (*aktu&#xFFFD; (*aktu&#xFFFD; (*aktu&#xFFFD; (*aktu&#xFFFD; (*aktu&#xFFFD; (*aktu&#xFFFD; (*aktu&#xFFFD; (*aktu&#xFFFD; (*aktu&#xFFFD; (*aktu&#xFFFD; (*aktu&#xFFFD; (*aktu&#xFFFD; (*aktu&#xFFFD; (*aktu&#xFFFD; (*aktu&#xFFFD; (*aktu&#xFFFD; (*aktu&#xFFFD; (*aktu&#xFFFD; (*aktu&#xFFFD; (*aktu&#xFFFD; (*aktu&#xFFFD; (*aktu&#xFFFD; (*aktu&#xFFFD; (*aktu&#xFFFD; (*aktu&#xFFFD; (*aktu&#xFFFD; (*aktu&#xFFFD; (*aktu&#xFFFD; (*aktu&#xFFFD; (*aktu&#xFFFD; (*aktu&#xFFFD; (*aktu&#xFFFD; (*aktu&#xFFFD; (*aktu&#xFFFD; (*aktu&#xFFFD; (*aktu&#xFFFD; (*aktu&#xFFFD; (*aktu&#xFFFD; (*aktu&#xFFFD; (*aktu&#xFFFD; (*aktu&#xFFFD; (*aktu&#xFFFD; (*aktu&#xFFFD; (*aktu&#xFFFD; (*aktu&#xFFFD; (*aktu&#xFFFD; (*aktu&#xFFFD; (*aktu&#xFFFD; (*aktu&#xFFFD; (*aktu&#xFFFD; (*aktu&#xFFFD; (*aktu&#xFFFD; (*aktu&#xFFFD; (*aktu&#xFFFD; (*aktu&#xFFFD; (*aktu&#xFFFD; (*aktu&#xFFFD; (*aktu&#xFFFD; (*aktu&#xFFFD; (*aktu&#xFFFD; (*aktu&#xFFFD; (*aktu&#xFFFD; (*aktu&#xFFFD; (*aktu&#xFFFD; (*aktu&#xFFFD; (*aktu&#xFFFD; (*aktu&#xFFFD; (*aktu&#xFFFD; (*aktu&#xFFFD; (*aktu&#xFFFD; (*aktu&#xFFFD; (*aktu&#xFFFD; (*aktu&#xFFFD; (*aktu&#xFFFD; (*aktu&#xFFFD; (*aktu&#xFFFD; (*aktu&#xFFFD; (*aktu&#xFFFD; (*aktu&#xFFFD; (*aktu&#xFFFD; (*aktu&#xFFFD; (*aktu&#xFFFD; (*aktu&#xFFFD; (*aktu&#xFFFD; (*aktu&#xFFFD; (*aktu&#xFFFD; (*aktu&#xFFFD; (*aktu&#xFFFD; (*aktu&#xFFFD; (*aktu&#xFFFD; (*aktu&#xFFFD; (*aktu&#xFFFD; (*aktu&#xFFFD; (*aktu&#xFFFD; (*aktu&#xFFFD; (*aktu&#xFFFD; (*aktu&#xFFFD; (*aktu&#xFFFD; (*aktu&#xFFFD; (*aktu&#xFFFD; (*aktu&#xFFFD; (*aktu&#xFFFD; (*aktu&#xFFFD; (*aktu&#xFFFD; (*aktu&#xFFFD; (*aktu&#xFFFD; (*aktu&#xFFFD; (*aktu&#xFFFD; (*aktu&#xFFFD; (*aktu&#xFFFD; (*aktu&#xFFFD; (*aktu&#xFFFD; (*aktu&#xFFFD; (*aktu&#xFFFD; (*aktu&#xFFFD; (*aktu&#xFFFD; (*aktu&#xFFFD; (*aktu&#xFFFD; (*aktu&#xFFFD; (*aktu&#xFFFD; (*aktu&#xFFFD; (*aktu&#xFFFD; (*aktu&#xFFFD; (*aktu&#xFFFD; (*aktu&#xFFFD; (*aktu&#xFFFD; (*aktu&#xFFFD; (*aktu&#xFFFD; (*aktu&#xFFFD; (*aktu&#xFFFD; (*aktu&#xFFFD; (*aktu&#xFFFD; (*aktu&#xFFFD; (*aktu&#xFFFD; (*aktu&#xFFFD; (*aktu&#xFFFD; (*aktu&#xFFFD; (*aktu&#xFFFD; (*aktu&#xFFFD; (*aktu&#xFFFD; (*aktu&#xFFFD; (*aktu&#xFFFD; (*aktu&#xFFFD; (*aktu&#xFFFD; (*aktu&#xFFFD; (*aktu&#xFFFD; (*aktu&#xFFFD; (*aktu&#xFFFD; (*aktu&#xFFFD; (*aktu&#xFFFD; (*aktu&#xFFFD; (*aktu&#xFFFD; (*aktu&#xFFFD; (*aktu&#xFFFD; (*aktu&#xFFFD; (*aktu&#xFFFD; (*aktu&#xFFFD; (*aktu&#xFFFD; (*aktu&#xFFFD; (*aktu&#xFFFD; (*aktu&#xFFFD; (*aktu&#xFFFD; (*aktu&#xFFFD; (*aktu&#xFFFD; (*aktu&#xFFFD; (*aktu&#xFFFD; (*aktu&#xFFFD; (*aktu&#xFFFD; (*aktu&#xFFFD; (*aktu&#xFFFD; (*aktu&#xFFFD; (*aktu&#xFFFD; (*aktu&#xFFFD; (*aktu&#xFFFD; (*aktu&#xFFFD; (*aktu&#xFFFD; (*aktu&#xFFFD; (*aktu&#xFFFD; (*aktu&#xFFFD; (*aktu&#xFFFD; (*aktu&#xFFFD; (*aktu&#xFFFD; (*aktu&#xFFFD; (*aktu&#xFFFD; (*aktu&#xFFFD; (*aktu&#xFFFD; (*aktu&#xFFFD; (*aktu&#xFFFD; (*aktu&#xFFFD; (*aktu&#xFFFD; (*aktu&#xFFFD; (*aktu&#xFFFD; (*aktu&#xFFFD; (*aktu&#xFFFD; (*aktu&#xFFFD; (*aktu&#xFFFD; (*aktu&#xFFFD; (*aktu&#xFFFD; (*aktu&#xFFFD; (*aktu&#xFFFD; (*aktu&#xFFFD; (*aktu&#xFFFD; (*aktu&#xFFFD; (*aktu&#xFFFD; (*aktu&#xFFFD; (*aktu&#xFFFD; (*aktu&#xFFFD; (*aktu&#xFFFD; (*aktu&#xFFFD; (*aktu&#xFFFD; (*aktu&#xFFFD; (*aktu&#xFFFD; (*aktu&#xFFFD; (*aktu&#xFFFD; (*aktu&#xFFFD; (*aktu&#xFFFD; (*aktu&#xFFFD; (*aktu&#xFFFD; (*aktu&#xFFFD; (*aktu&#xFFFD; (*aktu&#xFFFD; (*aktu&#xFFFD; (*aktu&#xFFFD; (*aktu&#xFFFD; (*aktu&#xFFFD; (*aktu&#xFFFD; (*aktu&#xFFFD; (*aktu&#xFFFD; (*aktu&#xFFFD; (*aktu&#xFFFD; (*aktu&#xFFFD; (*aktu&#xFFFD; (*aktu&#xFFFD; (*aktu&#xFFFD; (*aktu&#xFFFD; (*aktu&#xFFFD; (*aktu&#xFFFD; (*aktu&#xFFFD; (*aktu&#xFFFD; (*aktu&#xFFFD; (*aktu&#xFFFD; (*aktu&#xFFFD; (*aktu&#xFFFD; (*aktu&#xFFFD; (*aktu&#xFFFD; (*aktu&#xFFFD; (*aktu&#xFFFD; (*aktu&#xFFFD; (*aktu&#xFFFD; (*aktu&#xFFFD; (*aktu&#xFFFD; (*aktu&#xFFFD; (*aktu&#xFFFD; (*aktu&#xFFFD; (*aktu&#xFFFD; (*aktu&#xFFFD; (*aktu&#xFFFD; (*aktu&#xFFFD; (*aktu&#xFFFD; (*aktu&#xFFFD; (*aktu&#xFFFD; (*aktu&#xFFFD; (*aktu&#xFFFD; (*aktu&#xFFFD; (*aktu&#xFFFD; (*aktu&#xFFFD; (*aktu&#xFFFD; (*aktu&#xFFFD; (*aktu&#xFFFD; (*aktu&#xFFFD; (*aktu&#xFFFD; (*aktu&#xFFFD; (*aktu&#xFFFD; (*aktu&#xFFFD; (*aktu&#xFFFD; (*aktu&#xFFFD; (*aktu&#xFFFD; (*aktu&#xFFFD; (*aktu&#xFFFD; (*aktu&#xFFFD; (*aktu&#xFFFD; (*aktu&#xFFFD; (*aktu&#xFFFD; (*aktu&#xFFFD; (*aktu&#xFFFD; (*aktu&#xFFFD; (*aktu&#xFFFD; (*aktu&#xFFFD; (*aktu&#xFFFD; (*aktu&#xFFFD; (*aktu&#xFFFD; (*aktu&#xFFFD; (*aktu&#xFFFD; (*aktu&#xFFFD; (*aktu&#xFFFD; (*aktu&#xFFFD; (*aktu&#xFFFD; (*aktu&#xFFFD; (*aktu&#xFFFD; (*aktu&#xFFFD; (*aktu&#xFFFD; (*aktu&#xFFFD; (*aktu&#xFFFD; (*aktu&#xFFFD; (*aktu&#xFFFD; (*aktu&#xFFFD; (*aktu&#xFFFD; (*aktu&#xFFFD; (*aktu&#xFFFD; (*aktu&#xFFFD; (*aktu&#xFFFD; (*aktu&#xFFFD; (*aktu&#xFFFD; (*aktu&#xFFFD; (*aktu&#xFFFD; (*aktu&#xFFFD; (*aktu&#xFFFD; (*aktu&#xFFFD; (*aktu&#xFFFD; (*aktu&#xFFFD; (*aktu&#xFFFD; (*aktu&#xFFFD; (*aktu&#xFFFD; (*aktu&#xFFFD; (*aktu&#xFFFD; (*aktu&#xFFFD; (*aktu&#xFFFD; (*aktu&#xFFFD; (*aktu&#xFFFD; (*aktu&#xFFFD; (*aktu&#xFFFD; (*aktu&#xFFFD; (*aktu&#xFFFD; (*aktu&#xFFFD; (*aktu&#xFFFD; (*aktu&#xFFFD; (*aktu&#xFFFD; (*aktu&#xFFFD; (*aktu&#xFFFD; (*aktu&#xFFFD; (*aktu&#xFFFD; (*aktu&#xFFFD; (*aktu&#xFFFD; (*aktu&#xFFFD; (*aktu&#xFFFD; (*aktu&#xFFFD; (*aktu&#xFFFD; (*aktu&#xFFFD; (*aktu&#xFFFD; (*aktu&#xFFFD; (*aktu&#xFFFD; (*aktu&#xFFFD; (*aktu&#xFFFD; (*aktu&#xFFFD; (*aktu&#xFFFD; (*aktu&#xFFFD; (*aktu&#xFFFD; (*aktu&#xFFFD; (*aktu&#xFFFD; (*aktu&#xFFFD; (*aktu&#xFFFD; (*aktu&#xFFFD; (*aktu&#xFFFD; (*aktu&#xFFFD; (*aktu&#xFFFD; (*aktu&#xFFFD; (*aktu&#xFFFD; (*aktu&#xFFFD; (*aktu&#xFFFD; (*aktu&#xFFFD; (*aktu&#xFFFD; (*aktu&#xFFFD; (*aktu&#xFFFD; (*aktu&#xFFFD; (*aktu&#xFFFD; (*aktu&#xFFFD; (*aktu&#xFFFD; (*aktu&#xFFFD; (*aktu&#xFFFD; (*aktu&#xFFFD; (*aktu&#xFFFD; (*aktu&#xFFFD; (*aktu&#xFFFD; (*aktu&#xFFFD; (*aktu&#xFFFD; (*aktu&#xFFFD; (*aktu&#xFFFD; (*aktu&#xFFFD; (*aktu&#xFFFD; (*aktu&#xFFFD; (*aktu&#xFFFD; (*aktu&#xFFFD; (*aktu&#xFFFD; (*aktu&#xFFFD; (*aktu&#xFFFD; (*aktu&#xFFFD; (*aktu&#xFFFD; (*aktu&#xFFFD; (*aktu&#xFFFD; (*aktu&#xFFFD; (*aktu&#xFFFD; (*aktu&#xFFFD; (*aktu&#xFFFD; (*aktu&#xFFFD; (*aktu&#xFFFD; (*aktu&#xFFFD; (*aktu&#xFFFD; (*aktu&#xFFFD; (*aktu&#xFFFD; (*aktu&#xFFFD; (*aktu&#xFFFD; (*aktu&#xFFFD; (*aktu&#xFFFD; (*aktu&#xFFFD; (*aktu&#xFFFD; (*aktu&#xFFFD; (*aktu&#xFFFD; (*aktu&#xFFFD; (*aktu&#xFFFD; (*aktu&#xFFFD; (*aktu&#xFFFD; (*aktu&#xFFFD; (*aktu&#xFFFD; (*aktu&#xFFFD; (*aktu&#xFFFD; (*aktu&#xFFFD; (*aktu&#xFFFD; (*aktu&#xFFFD; (*aktu&#xFFFD; (*aktu&#xFFFD; (*aktu&#xFFFD; (*aktu&#xFFFD; (*aktu&#xFFFD; (*aktu&#xFFFD; (*aktu&#xFFFD; (*aktu&#xFFFD; (*aktu&#xFFFD; (*aktu&#xFFFD; (*aktu&#xFFFD; (*aktu&#xFFFD; (*aktu&#xFFFD; (*aktu&#xFFFD; (*aktu&#xFFFD; (*aktu&#xFFFD; (*aktu&#xFFFD; (*aktu&#xFFFD; (*aktu&#xFFFD; (*aktu&#xFFFD; (*aktu&#xFFFD; (*aktu&#xFFFD; (*aktu&#xFFFD; (*aktu&#xFFFD; (*aktu&#xFFFD; (*aktu&#xFFFD; (*aktu&#xFFFD; (*aktu&#xFFFD; (*aktu&#xFFFD; (*aktu&#xFFFD; (*aktu&#xFFFD; (*aktu&#xFFFD; (*aktu&#xFFFD; (*aktu&#xFFFD; (*aktu&#xFFFD; (*aktu&#xFFFD; (*aktu&#xFFFD; (*aktu&#xFFFD; (*aktu&#xFFFD; (*aktu&#xFFFD; (*aktu&#xFFFD; (*aktu&#xFFFD; (*aktu&#xFFFD; (*aktu&#xFFFD; (*aktu&#xFFFD; (*aktu&#xFFFD; (*aktu&#xFFFD; (*aktu&#xFFFD; (*aktu&#xFFFD; (*aktu&#xFFFD; (*aktu&#xFFFD; (*aktu&#xFFFD; (*aktu&#xFFFD; (*aktu&#xFFFD; (*aktu&#xFFFD; (*aktu&#xFFFD; (*aktu&#xFFFD; (*aktu&#xFFFD; (*aktu&#xFFFD; (*aktu&#xFFFD; (*aktu&#xFFFD; (*aktu&#xFFFD; (*aktu&#xFFFD; (*aktu&#xFFFD; (*aktu&#xFFFD; (*aktu&#xFFFD; (*aktu&#xFFFD; (*aktu&#xFFFD; (*aktu&#xFFFD; (*aktu&#xFFFD; (*aktu&#xFFFD; (*aktu&#xFFFD; (*aktu&#xFFFD; (*aktu&#xFFFD; (*aktu&#xFFFD; (*aktu&#xFFFD; (*aktu&#xFFFD; (*aktu&#xFFFD; (*aktu&#xFFFD; (*aktu&#xFFFD; (*aktu&#xFFFD; (*aktu&#xFFFD; (*aktu&#xFFFD; (*aktu&#xFFFD; (*aktu&#xFFFD; (*aktu&#xFFFD; (*aktu&#xFFFD; (*aktu&#xFFFD; (*aktu&#xFFFD; (*aktu&#xFFFD; (*aktu&#xFFFD; (*aktu&#xFFFD; (*aktu&#xFFFD; (*aktu&#xFFFD; (*aktu&#xFFFD; (*aktu&#xFFFD; (*aktu&#xFFFD; (*aktu&#xFFFD; (*aktu&#xFFFD; (*aktu&#xFFFD; (*aktu&#xFFFD; (*aktu&#xFFFD; (*aktu&#xFFFD; (*aktu&#xFFFD; (*aktu&#xFFFD; (*aktu&#xFFFD; (*aktu&#xFFFD; (*aktu&#xFFFD; (*aktu&#xFFFD; (*aktu&#xFFFD; (*aktu&#xFFFD; (*aktu&#xFFFD; (*aktu&#xFFFD; (*aktu&#xFFFD; (*aktu&#xFFFD; (*aktu&#xFFFD; (*aktu&#xFFFD; (*aktu&#xFFFD; (*aktu&#xFFFD; (*aktu&#xFFFD; (*aktu&#xFFFD; (*aktu&#xFFFD; (*aktu&#xFFFD; (*aktu&#xFFFD; (*aktu&#xFFFD; (*aktu&#xFFFD; (*aktu&#xFFFD; (*aktu&#xFFFD; (*aktu&#xFFFD; (*aktu&#xFFFD; (*aktu&#xFFFD; (*aktu&#xFFFD; (*aktu&#xFFFD; (*aktu&#xFFFD; (*aktu&#xFFFD; (*aktu&#xFFFD; (*aktu&#xFFFD; (*aktu&#xFFFD; (*aktu&#xFFFD; (*aktu&#xFFFD; (*aktu&#xFFFD; (*aktu&#xFFFD; (*aktu&#xFFFD; (*aktu&#xFFFD; (*aktu&#xFFFD; (*aktu&#xFFFD; (*aktu&#xFFFD; (*aktu&#xFFFD; (*aktu&#xFFFD; (*aktu&#xFFFD; (*aktu&#xFFFD; (*aktu&#xFFFD; (*aktu&#xFFFD; (*aktu&#xFFFD; (*aktu&#xFFFD; (*aktu&#xFFFD; (*aktu&#xFFFD; (*aktu&#xFFFD; (*aktu&#xFFFD; (*aktu&#xFFFD; (*aktu&#xFFFD; (*aktu&#xFFFD; (*aktu&#xFFFD; (*aktu&#xFFFD; (*aktu&#xFFFD; (*aktu&#xFFFD; (*aktu&#xFFFD; (*aktu&#xFFFD; (*aktu&#xFFFD; (*aktu&#xFFFD; (*aktu&#xFFFD; (*aktu&#xFFFD; (*aktu&#xFFFD; (*aktu&#xFFFD; (*aktu&#xFFFD; (*aktu&#xFFFD; (*aktu&#xFFFD; (*aktu&#xFFFD; (*aktu&#xFFFD; (*aktu&#xFFFD; (*aktu&#xFFFD; (*aktu&#xFFFD; (*aktu&#xFFFD; (*aktu&#xFFFD; (*aktu&#xFFFD; (*aktu&#xFFFD; (*aktu&#xFFFD; (*aktu&#xFFFD; (*aktu&#xFFFD; (*aktu&#xFFFD; (*aktu&#xFFFD; (*aktu&#xFFFD; (*aktu&#xFFFD; (*aktu&#xFFFD; (*aktu&#xFFFD; (*aktu&#xFFFD; (*aktu&#xFFFD; (*aktu&#xFFFD; (*aktu&#xFFFD; (*aktu&#xFFFD; (*aktu&#xFFFD; (*aktu&#xFFFD; (*aktu&#xFFFD; (*aktu&#xFFFD; (*aktu&#xFFFD; (*aktu&#xFFFD; (*aktu&#xFFFD; (*aktu&#xFFFD; (*aktu&#xFFFD; (*aktu&#xFFFD; (*aktu&#xFFFD; (*aktu&#xFFFD; (*aktu&#xFFFD; (*aktu&#xFFFD; (*aktu&#xFFFD; (*aktu&#xFFFD; (*aktu&#xFFFD; (*aktu&#xFFFD; (*aktu&#xFFFD; (*aktu&#xFFFD; (*aktu&#xFFFD; (*aktu&#xFFFD; (*aktu&#xFFFD; (*aktu&#xFFFD; (*aktu&#xFFFD; (*aktu&#xFFFD; (*aktu&#xFFFD; (*aktu&#xFFFD; (*aktu&#xFFFD; (*aktu&#xFFFD; (*aktu&#xFFFD; (*aktu&#xFFFD; (*aktu&#xFFFD; (*aktu&#xFFFD; (*aktu&#xFFFD; (*aktu&#xFFFD; (*aktu&#xFFFD; (*aktu&#xFFFD; (*aktu&#xFFFD; (*aktu&#xFFFD; (*aktu&#xFFFD; (*aktu&#xFFFD; (*aktu&#xFFFD; (*aktu&#xFFFD; (*aktu&#xFFFD; (*aktu&#xFFFD; (*aktu&#xFFFD; (*aktu&#xFFFD; (*aktu&#xFFFD; (*aktu&#xFFFD; (*aktu&#xFFFD; (*aktu&#xFFFD; (*aktu&#xFFFD; (*aktu&#xFFFD; (*aktu&#xFFFD; (*aktu&#xFFFD; (*aktu&#xFFFD; (*aktu&#xFFFD; (*aktu&#xFFFD; (*aktu&#xFFFD; (*aktu&#xFFFD; (*aktu&#xFFFD; (*aktu&#xFFFD; (*aktu&#xFFFD; (*aktu&#xFFFD; (*aktu&#xFFFD; (*aktu&#xFFFD; (*aktu&#xFFFD; (*aktu&#xFFFD; (*aktu&#xFFFD; (*aktu&#xFFFD; (*aktu&#xFFFD; (*aktu&#xFFFD; (*aktu&#xFFFD; (*aktu&#xFFFD; (*aktu&#xFFFD; (*aktu&#xFFFD; (*aktu&#xFFFD; (*aktu&#xFFFD; (*aktu&#xFFFD; (*aktu&#xFFFD; (*aktu&#xFFFD; (*aktu&#xFFFD; (*aktu&#xFFFD; (*aktu&#xFFFD; (*aktu&#xFFFD; (*aktu&#xFFFD; (*aktu&#xFFFD; (*aktu&#xFFFD; (*aktu&#xFFFD; (*aktu&#xFFFD; (*aktu&#xFFFD; (*aktu&#xFFFD; (*aktu&#xFFFD; (*aktu&#xFFFD; (*aktu&#xFFFD; (*aktu&#xFFFD; (*aktu&#xFFFD; (*aktu&#xFFFD; (*aktu&#xFFFD; (*aktu&#xFFFD; (*aktu&#xFFFD; (*aktu&#xFFFD; (*aktu&#xFFFD; (*aktu&#xFFFD; (*aktu&#xFFFD; (*aktu&#xFFFD; (*aktu&#xFFFD; (*aktu&#xFFFD; (*aktu&#xFFFD; (*aktu&#xFFFD; (*aktu&#xFFFD; (*aktu&#xFFFD; (*aktu&#xFFFD; (*aktu&#xFFFD; (*aktu&#xFFFD; (*aktu&#xFFFD; (*aktu&#xFFFD; (*aktu&#xFFFD; (*aktu&#xFFFD; (*aktu&#xFFFD; (*aktu&#xFFFD; (*aktu&#xFFFD; (*aktu&#xFFFD; (*aktu&#xFFFD; (*aktu&#xFFFD; (*aktu&#xFFFD; (*aktu&#xFFFD; (*aktu&#xFFFD; (*aktu&#xFFFD; (*aktu&#xFFFD; (*aktu&#xFFFD; (*aktu&#xFFFD; (*aktu&#xFFFD; (*aktu&#xFFFD; (*aktu&#xFFFD; (*aktu&#xFFFD; (*aktu&#xFFFD; (*aktu&#xFFFD; (*aktu&#xFFFD; (*aktu&#xFFFD; (*aktu&#xFFFD; (*aktu&#xFFFD; (*aktu&#xFFFD; (*aktu&#xFFFD; (*aktu&#xFFFD; (*aktu&#xFFFD; (*aktu&#xFFFD; (*aktu&#xFFFD; (*aktu&#xFFFD; (*aktu&#xFFFD; (*aktu&#xFFFD; (*aktu&#xFFFD; (*aktu&#xFFFD; (*aktu&#xFFFD; (*aktu&#xFFFD; (*aktu&#xFFFD; (*aktu&#xFFFD; (*aktu&#xFFFD; (*aktu&#xFFFD; (*aktu&#xFFFD; (*aktu&#xFFFD; (*aktu&#xFFFD; (*aktu&#xFFFD; (*aktu&#xFFFD; (*aktu&#xFFFD; (*aktu&#xFFFD; (*aktu&#xFFFD; (*aktu&#xFFFD; (*aktu&#xFFFD; (*aktu&#xFFFD; (*aktu&#xFFFD; (*aktu&#xFFFD; (*aktu&#xFFFD; (*aktu&#xFFFD; (*aktu&#xFFFD; (*aktu&#xFFFD; (*aktu&#xFFFD; (*aktu&#xFFFD; (*aktu&#xFFFD; (*aktu&#xFFFD; (*aktu&#xFFFD; (*aktu&#xFFFD; (*aktu&#xFFFD; (*aktu&#xFFFD; (*aktu&#xFFFD; (*aktu&#xFFFD; (*aktu&#xFFFD; (*aktu&#xFFFD; (*aktu&#xFFFD; (*aktu&#xFFFD; (*aktu&#xFFFD; (*aktu&#xFFFD; (*aktu&#xFFFD; (*aktu&#xFFFD; (*aktu&#xFFFD; (*aktu&#xFFFD; (*aktu&#xFFFD; (*aktu&#xFFFD; (*aktu&#xFFFD; (*aktu&#xFFFD; (*aktu&#xFFFD; (*aktu&#xFFFD; (*aktu&#xFFFD; (*aktu&#xFFFD; (*aktu&#xFFFD; (*aktu&#xFFFD; (*aktu&#xFFFD; (*aktu&#xFFFD; (*aktu&#xFFFD; (*aktu&#xFFFD; (*aktu&#xFFFD; (*aktu&#xFFFD; (*aktu&#xFFFD; (*aktu&#xFFFD; (*aktu&#xFFFD; (*aktu&#xFFFD; (*aktu&#xFFFD; (*aktu&#xFFFD; (*aktu&#xFFFD; (*aktu&#xFFFD; (*aktu&#xFFFD; (*aktu&#xFFFD; (*aktu&#xFFFD; (*aktu&#xFFFD; (*aktu&#xFFFD; (*aktu&#xFFFD; (*aktu&#xFFFD; (*aktu&#xFFFD; (*aktu&#xFFFD; (*aktu&#xFFFD; (*aktu&#xFFFD; (*aktu&#xFFFD; (*aktu&#xFFFD; (*aktu&#xFFFD; (*aktu&#xFFFD; (*aktu&#xFFFD; (*aktu&#xFFFD; (*aktu&#xFFFD; (*aktu&#xFFFD; (*aktu&#xFFFD; (*aktu&#xFFFD; (*aktu&#xFFFD; (*aktu&#xFFFD; (*aktu&#xFFFD; (*aktu&#xFFFD; (*aktu&#xFFFD; (*aktu&#xFFFD; (*aktu&#xFFFD; (*aktu&#xFFFD; (*aktu&#xFFFD; (*aktu&#xFFFD; (*aktu&#xFFFD; (*aktu&#xFFFD; (*aktu&#xFFFD; (*aktu&#xFFFD; (*aktu&#xFFFD; (*aktu&#xFFFD; (*aktu&#xFFFD; (*aktu&#xFFFD; (*aktu&#xFFFD; (*aktu&#xFFFD; (*aktu&#xFFFD; (*aktu&#xFFFD; (*aktu&#xFFFD; (*aktu&#xFFFD; (*aktu&#xFFFD; (*aktu&#xFFFD; (*aktu&#xFFFD; (*aktu&#xFFFD; (*aktu&#xFFFD; (*aktu&#xFFFD; (*aktu&#xFFFD; (*aktu&#xFFFD; (*aktu&#xFFFD; (*aktu&#xFFFD; (*aktu&#xFFFD; (*aktu&#xFFFD; (*aktu&#xFFFD; (*aktu&#xFFFD; (*aktu&#xFFFD; (*aktu&#xFFFD; (*aktu&#xFFFD; (*aktu&#xFFFD; (*aktu&#xFFFD; (*aktu&#xFFFD; (*aktu&#xFFFD; (*aktu&#xFFFD; (*aktu&#xFFFD; (*aktu&#xFFFD; (*aktu&#xFFFD; (*aktu&#xFFFD; (*aktu&#xFFFD; (*aktu&#xFFFD; (*aktu&#xFFFD; (*aktu&#xFFFD; (*aktu&#xFFFD; (*aktu&#xFFFD; (*aktu&#xFFFD; (*aktu&#xFFFD; (*aktu&#xFFFD; (*aktu&#xFFFD; (*aktu&#xFFFD; (*aktu&#xFFFD; (*aktu&#xFFFD; (*aktu&#xFFFD; (*aktu&#xFFFD; (*aktu&#xFFFD; (*aktu&#xFFFD; (*aktu&#xFFFD; (*aktu&#xFFFD; (*aktu&#xFFFD; (*aktu&#xFFFD; (*aktu&#xFFFD; (*aktu&#xFFFD; (*aktu&#xFFFD; (*aktu&#xFFFD; (*aktu&#xFFFD; (*aktu&#xFFFD; (*aktu&#xFFFD; (*aktu&#xFFFD; (*aktu&#xFFFD; (*aktu&#xFFFD; (*aktu&#xFFFD; (*aktu&#xFFFD; (*aktu&#xFFFD; (*aktu&#xFFFD; (*aktu&#xFFFD; (*aktu&#xFFFD; (*aktu&#xFFFD; (*aktu&#xFFFD; (*aktu&#xFFFD; (*aktu&#xFFFD; (*aktu&#xFFFD; (*aktu&#xFFFD; (*aktu&#xFFFD; (*aktu&#xFFFD; (*aktu&#xFFFD; (*aktu&#xFFFD; (*aktu&#xFFFD; (*aktu&#xFFFD; (*aktu&#xFFFD; (*aktu&#xFFFD; (*aktu&#xFFFD; (*aktu&#xFFFD; (*aktu&#xFFFD; (*aktu&#xFFFD; (*aktu&#xFFFD; (*aktu&#xFFFD; (*aktu&#xFFFD; (*aktu&#xFFFD; (*aktu&#xFFFD; (*aktu&#xFFFD; (*aktu&#xFFFD; (*aktu&#xFFFD; (*aktu&#xFFFD; (*aktu&#xFFFD; (*aktu&#xFFFD; (*aktu&#xFFFD; (*aktu&#xFFFD; (*aktu&#xFFFD; (*aktu&#xFFFD; (*aktu&#xFFFD; (*aktu&#xFFFD; (*aktu&#xFFFD; (*aktu&#xFFFD; (*aktu&#xFFFD; (*aktu&#xFFFD; (*aktu&#xFFFD; (*aktu&#xFFFD; (*aktu&#xFFFD; (*aktu&#xFFFD; (*aktu&#xFFFD; (*aktu&#xFFFD; (*aktu&#xFFFD; (*aktu&#xFFFD; (*aktu&#xFFFD; (*aktu&#xFFFD; (*aktu&#xFFFD; (*aktu&#xFFFD; (*aktu&#xFFFD; (*aktu&#xFFFD; (*aktu&#xFFFD; (*aktu&#xFFFD; (*aktu&#xFFFD; (*aktu&#xFFFD; (*aktu&#xFFFD; (*aktu&#xFFFD; (*aktu&#xFFFD; (*aktu&#xFFFD; (*aktu&#xFFFD; (*aktu&#xFFFD; (*aktu&#xFFFD; (*aktu&#xFFFD; (*aktu&#xFFFD; (*aktu&#xFFFD; (*aktu&#xFFFD; (*aktu&#xFFFD; (*aktu&#xFFFD; (*aktu&#xFFFD; (*aktu&#xFFFD; (*aktu&#xFFFD; (*aktu&#xFFFD; (*aktu&#xFFFD; (*aktu&#xFFFD; (*aktu&#xFFFD; (*aktu&#xFFFD; (*aktu&#xFFFD; (*aktu&#xFFFD; (*aktu&#xFFFD; (*aktu&#xFFFD; (*aktu&#xFFFD; (*aktu&#xFFFD; (*aktu&#xFFFD; (*aktu&#xFFFD; (*aktu&#xFFFD; (*aktu&#xFFFD; (*aktu&#xFFFD; (*aktu&#xFFFD; (*aktu&#xFFFD; (*aktu&#xFFFD; (*aktu&#xFFFD; (*aktu&#xFFFD; (*aktu&#xFFFD; (*aktu&#xFFFD; (*aktu&#xFFFD; (*aktu&#xFFFD; (*aktu&#xFFFD; (*aktu&#xFFFD; (*aktu&#xFFFD; (*aktu&#xFFFD; (*aktu&#xFFFD; (*aktu&#xFFFD; (*aktu&#xFFFD; (*aktu&#xFFFD; (*aktu&#xFFFD; (*aktu&#xFFFD; (*aktu&#xFFFD; (*aktu&#xFFFD; (*aktu&#xFFFD; (*aktu&#xFFFD; (*aktu&#xFFFD; (*aktu&#xFFFD; (*aktu&#xFFFD; (*aktu&#xFFFD; (*aktu&#xFFFD; (*aktu&#xFFFD; (*aktu&#xFFFD; (*aktu&#xFFFD; (*aktu&#xFFFD; (*aktu&#xFFFD; (*aktu&#xFFFD; (*aktu&#xFFFD; (*aktu&#xFFFD; (*aktu&#xFFFD; (*aktu&#xFFFD; (*aktu&#xFFFD; (*aktu&#xFFFD; (*aktu&#xFFFD; (*aktu&#xFFFD; (*aktu&#xFFFD; (*aktu&#xFFFD; (*aktu&#xFFFD; (*aktu&#xFFFD; (*aktu&#xFFFD; (*aktu&#xFFFD; (*aktu&#xFFFD; (*aktu&#xFFFD; (*aktu&#xFFFD; (*aktu&#xFFFD; (*aktu&#xFFFD; (*aktu&#xFFFD; (*aktu&#xFFFD; (*aktu&#xFFFD; (*aktu&#xFFFD; (*aktu&#xFFFD; (*aktu&#xFFFD; (*aktu&#xFFFD; (*aktu&#xFFFD; (*aktu&#xFFFD; (*aktu&#xFFFD; (*aktu&#xFFFD; (*aktu&#xFFFD; (*aktu&#xFFFD; (*aktu&#xFFFD; (*aktu&#xFFFD; (*aktu&#xFFFD; (*aktu&#xFFFD; (*aktu&#xFFFD; (*aktu&#xFFFD; (*aktu&#xFFFD; (*aktu&#xFFFD; (*aktu&#xFFFD; (*aktu&#xFFFD; (*aktu&#xFFFD; (*aktu&#xFFFD; (*aktu&#xFFFD; (*aktu&#xFFFD; (*aktu&#xFFFD; (*aktu&#xFFFD; (*aktu&#xFFFD; (*aktu&#xFFFD; (*aktu&#xFFFD; (*aktu&#xFFFD; (*aktu&#xFFFD; (*aktu&#xFFFD; (*aktu&#xFFFD; (*aktu&#xFFFD; (*aktu&#xFFFD; (*aktu&#xFFFD; (*aktu&#xFFFD; (*aktu&#xFFFD; (*aktu&#xFFFD; (*aktu&#xFFFD; (*aktu&#xFFFD; (*aktu&#xFFFD; (*aktu&#xFFFD; (*aktu&#xFFFD; (*aktu&#xFFFD; (*aktu&#xFFFD; (*aktu&#xFFFD; (*aktu&#xFFFD; (*aktu&#xFFFD; (*aktu&#xFFFD; (*aktu&#xFFFD; (*aktu&#xFFFD; (*aktu&#xFFFD; (*aktu&#xFFFD; (*aktu&#xFFFD; (*aktu&#xFFFD; (*aktu&#xFFFD; (*aktu&#xFFFD; (*aktu&#xFFFD; (*aktu&#xFFFD; (*aktu&#xFFFD; (*aktu&#xFFFD; (*aktu&#xFFFD; (*aktu&#xFFFD; (*aktu&#xFFFD; (*aktu&#xFFFD; (*aktu&#xFFFD; (*aktu&#xFFFD; (*aktu&#xFFFD; (*aktu&#xFFFD; (*aktu&#xFFFD; (*aktu&#xFFFD; (*aktu&#xFFFD; (*aktu&#xFFFD; (*aktu&#xFFFD; (*aktu&#xFFFD; (*aktu&#xFFFD; (*aktu&#xFFFD; (*aktu&#xFFFD; (*aktu&#xFFFD; (*aktu&#xFFFD; (*aktu&#xFFFD; (*aktu&#xFFFD; (*aktu&#xFFFD; (*aktu&#xFFFD; (*aktu&#xFFFD; (*aktu&#xFFFD; (*aktu&#xFFFD; (*aktu&#xFFFD; (*aktu&#xFFFD; (*aktu&#xFFFD; (*aktu&#xFFFD; (*aktu&#xFFFD; (*aktu&#xFFFD; (*aktu&#xFFFD; (*aktu&#xFFFD; (*aktu&#xFFFD; (*aktu&#xFFFD; (*aktu&#xFFFD; (*aktu&#xFFFD; (*aktu&#xFFFD; (*aktu&#xFFFD; (*aktu&#xFFFD; (*aktu&#xFFFD; (*aktu&#xFFFD; (*aktu&#xFFFD; (*aktu&#xFFFD; (*aktu&#xFFFD; (*aktu&#xFFFD; (*aktu&#xFFFD; (*aktu&#xFFFD; (*aktu&#xFFFD; (*aktu&#xFFFD; (*aktu&#xFFFD; (*aktu&#xFFFD; (*aktu&#xFFFD; (*aktu&#xFFFD; (*aktu&#xFFFD; (*aktu&#xFFFD; (*aktu&#xFFFD; (*aktu&#xFFFD; (*aktu&#xFFFD; (*aktu&#xFFFD; (*aktu&#xFFFD; (*aktu&#xFFFD; (*aktu&#xFFFD; (*aktu&#xFFFD; (*aktu&#xFFFD; (*aktu&#xFFFD; (*aktu&#xFFFD; (*aktu&#xFFFD; (*aktu&#xFFFD; (*aktu&#xFFFD; (*aktu&#xFFFD; (*aktu&#xFFFD; (*aktu&#xFFFD; (*aktu&#xFFFD; (*aktu&#xFFFD; (*aktu&#xFFFD; (*aktu&#xFFFD; (*aktu&#xFFFD; (*aktu&#xFFFD; (*aktu&#xFFFD; (*aktu&#xFFFD; (*aktu&#xFFFD; (*aktu&#xFFFD; (*aktu&#xFFFD; (*aktu&#xFFFD; (*aktu&#xFFFD; (*aktu&#xFFFD; (*aktu&#xFFFD; (*aktu&#xFFFD; (*aktu&#xFFFD; (*aktu&#xFFFD; (*aktu&#xFFFD; (*aktu&#xFFFD; (*aktu&#xFFFD; (*aktu&#xFFFD; (*aktu&#xFFFD; (*aktu&#xFFFD; (*aktu&#xFFFD; (*aktu&#xFFFD; (*aktu&#xFFFD; (*aktu&#xFFFD; (*aktu&#xFFFD; (*aktu&#xFFFD; (*aktu&#xFFFD; (*aktu&#xFFFD; (*aktu&#xFFFD; (*aktu&#xFFFD; (*aktu&#xFFFD; (*aktu&#xFFFD; (*aktu&#xFFFD; (*aktu&#xFFFD; (*aktu&#xFFFD; (*aktu&#xFFFD; (*aktu&#xFFFD; (*aktu&#xFFFD; (*aktu&#xFFFD; (*aktu&#xFFFD; (*aktu&#xFFFD; (*aktu&#xFFFD; (*aktu&#xFFFD; (*aktu&#xFFFD; (*aktu&#xFFFD; (*aktu&#xFFFD; (*aktu&#xFFFD; (*aktu&#xFFFD; (*aktu&#xFFFD; (*aktu&#xFFFD; (*aktu&#xFFFD; (*aktu&#xFFFD; (*aktu&#xFFFD; (*aktu&#xFFFD; (*aktu&#xFFFD; (*aktu&#xFFFD; (*aktu&#xFFFD; (*aktu&#xFFFD; (*aktu&#xFFFD; (*aktu&#xFFFD; (*aktu&#xFFFD; (*aktu&#xFFFD; (*aktu&#xFFFD; (*aktu&#xFFFD; (*aktu&#xFFFD; (*aktu&#xFFFD; (*aktu&#xFFFD; (*aktu&#xFFFD; (*aktu&#xFFFD; (*aktu&#xFFFD; (*aktu&#xFFFD; (*aktu&#xFFFD; (*aktu&#xFFFD; (*aktu&#xFFFD; (*aktu&#xFFFD; (*aktu&#xFFFD; (*aktu&#xFFFD; (*aktu&#xFFFD; (*aktu&#xFFFD; (*aktu&#xFFFD; (*aktu&#xFFFD; (*aktu&#xFFFD; (*aktu&#xFFFD; (*aktu&#xFFFD; (*aktu&#xFFFD; (*aktu&#xFFFD; (*aktu&#xFFFD; (*aktu&#xFFFD; (*aktu&#xFFFD; (*aktu&#xFFFD; (*aktu&#xFFFD; (*aktu&#xFFFD; (*aktu&#xFFFD; (*aktu&#xFFFD; (*aktu&#xFFFD; (*aktu&#xFFFD; (*aktu&#xFFFD; (*aktu&#xFFFD; (*aktu&#xFFFD; (*aktu&#xFFFD; (*aktu&#xFFFD; (*aktu&#xFFFD; (*aktu&#xFFFD; (*aktu&#xFFFD; (*aktu&#xFFFD; (*aktu&#xFFFD; (*aktu&#xFFFD; (*aktu&#xFFFD; (*aktu&#xFFFD; (*aktu&#xFFFD; (*aktu&#xFFFD; (*aktu&#xFFFD; (*aktu&#xFFFD; (*aktu&#xFFFD; (*aktu&#xFFFD; (*aktu&#xFFFD; (*aktu&#xFFFD; (*aktu&#xFFFD; (*aktu&#xFFFD; (*aktu&#xFFFD; (*aktu&#xFFFD; (*aktu&#xFFFD; (*aktu&#xFFFD; (*aktu&#xFFFD; (*aktu&#xFFFD; (*aktu&#xFFFD; (*aktu&#xFFFD; (*aktu&#xFFFD; (*aktu&#xFFFD; (*aktu&#xFFFD; (*aktu&#xFFFD; (*aktu&#xFFFD; (*aktu&#xFFFD; (*aktu&#xFFFD; (*aktu&#xFFFD; (*aktu&#xFFFD; (*aktu&#xFFFD; (*aktu&#xFFFD; (*aktu&#xFFFD; (*aktu&#xFFFD; (*aktu&#xFFFD; (*aktu&#xFFFD; (*aktu&#xFFFD; (*aktu&#xFFFD; (*aktu&#xFFFD; (*aktu&#xFFFD; (*aktu&#xFFFD; (*aktu&#xFFFD; (*aktu&#xFFFD; (*aktu&#xFFFD; (*aktu&#xFFFD; (*aktu&#xFFFD; (*aktu&#xFFFD; (*aktu&#xFFFD; (*aktu&#xFFFD; (*aktu&#xFFFD; (*aktu&#xFFFD; (*aktu&#xFFFD; (*aktu&#xFFFD; (*aktu&#xFFFD; (*aktu&#xFFFD; (*aktu&#xFFFD; (*aktu&#xFFFD; (*aktu&#xFFFD; (*aktu&#xFFFD; (*aktu&#xFFFD; (*aktu&#xFFFD; (*aktu&#xFFFD; (*aktu&#xFFFD; (*aktu&#xFFFD; (*aktu&#xFFFD; (*aktu&#xFFFD; (*aktu&#xFFFD; (*aktu&#xFFFD; (*aktu&#xFFFD; (*aktu&#xFFFD; (*aktu&#xFFFD; (*aktu&#xFFFD; (*aktu&#xFFFD; (*aktu&#xFFFD; (*aktu&#xFFFD; (*aktu&#xFFFD; (*aktu&#xFFFD; (*aktu&#xFFFD; (*aktu&#xFFFD; (*aktu&#xFFFD; (*aktu&#xFFFD; (*aktu&#xFFFD; (*aktu&#xFFFD; (*aktu&#xFFFD; (*aktu&#xFFFD; (*aktu&#xFFFD; (*aktu&#xFFFD; (*aktu&#xFFFD; (*aktu&#xFFFD; (*aktu&#xFFFD; (*aktu&#xFFFD; (*aktu&#xFFFD; (*aktu&#xFFFD; (*aktu&#xFFFD; (*aktu&#xFFFD; (*aktu&#xFFFD; (*aktu&#xFFFD; (*aktu&#xFFFD; (*aktu&#xFFFD; (*aktu&#xFFFD; (*aktu&#xFFFD; (*aktu&#xFFFD; (*aktu&#xFFFD; (*aktu&#xFFFD; (*aktu&#xFFFD; (*aktu&#xFFFD; (*aktu&#xFFFD; (*aktu&#xFFFD; (*aktu&#xFFFD; (*aktu&#xFFFD; (*aktu&#xFFFD; (*aktu&#xFFFD; (*aktu&#xFFFD; (*aktu&#xFFFD; (*aktu&#xFFFD; (*aktu&#xFFFD; (*aktu&#xFFFD; (*aktu&#xFFFD; (*aktu&#xFFFD; (*aktu&#xFFFD; (*aktu&#xFFFD; (*aktu&#xFFFD; (*aktu&#xFFFD; (*aktu&#xFFFD; (*aktu&#xFFFD; (*aktu&#xFFFD; (*aktu&#xFFFD; (*aktu&#xFFFD; (*aktu&#xFFFD; (*aktu&#xFFFD; (*aktu&#xFFFD; (*aktu&#xFFFD; (*aktu&#xFFFD; (*aktu&#xFFFD; (*aktu&#xFFFD; (*aktu&#xFFFD; (*aktu&#xFFFD; (*aktu&#xFFFD; (*aktu&#xFFFD; (*aktu&#xFFFD; (*aktu&#xFFFD; (*aktu&#xFFFD; (*aktu&#xFFFD; (*aktu&#xFFFD; (*aktu&#xFFFD; (*aktu&#xFFFD; (*aktu&#xFFFD; (*aktu&#xFFFD; (*aktu&#xFFFD; (*aktu&#xFFFD; (*aktu&#xFFFD; (*aktu&#xFFFD; (*aktu&#xFFFD; (*aktu&#xFFFD; (*aktu&#xFFFD; (*aktu&#xFFFD; (*aktu&#xFFFD; (*aktu&#xFFFD; (*aktu&#xFFFD; (*aktu&#xFFFD; (*aktu&#xFFFD; (*aktu&#xFFFD; (*aktu&#xFFFD; (*aktu&#xFFFD; (*aktu&#xFFFD; (*aktu&#xFFFD; (*aktu&#xFFFD; (*aktu&#xFFFD; (*aktu&#xFFFD; (*aktu&#xFFFD; (*aktu&#xFFFD; (*aktu&#xFFFD; (*aktu&#xFFFD; (*aktu&#xFFFD; (*aktu&#xFFFD; (*aktu&#xFFFD; (*aktu&#xFFFD; (*aktu&#xFFFD; (*aktu&#xFFFD; (*aktu&#xFFFD; (*aktu&#xFFFD; (*aktu&#xFFFD; (*aktu&#xFFFD; (*aktu&#xFFFD; (*aktu&#xFFFD; (*aktu&#xFFFD; (*aktu&#xFFFD; (*aktu&#xFFFD; (*aktu&#xFFFD; (*aktu&#xFFFD; (*aktu&#xFFFD; (*aktu&#xFFFD; (*aktu&#xFFFD; (*aktu&#xFFFD; (*aktu&#xFFFD; (*aktu&#xFFFD; (*aktu&#xFFFD; (*aktu&#xFFFD; (*aktu&#xFFFD; (*aktu&#xFFFD; (*aktu&#xFFFD; (*aktu&#xFFFD; (*aktu&#xFFFD; (*aktu&#xFFFD; (*aktu&#xFFFD; (*aktu&#xFFFD; (*aktu&#xFFFD; (*aktu&#xFFFD; (*aktu&#xFFFD; (*aktu&#xFFFD; (*aktu&#xFFFD; (*aktu&#xFFFD; (*aktu&#xFFFD; (*aktu&#xFFFD; (*aktu&#xFFFD; (*aktu&#xFFFD; (*aktu&#xFFFD; (*aktu&#xFFFD; (*aktu&#xFFFD; (*aktu&#xFFFD; (*aktu&#xFFFD; (*aktu&#xFFFD; (*aktu&#xFFFD; (*aktu&#xFFFD; (*aktu&#xFFFD; (*aktu&#xFFFD; (*aktu&#xFFFD; (*aktu&#xFFFD; (*aktu&#xFFFD; (*aktu&#xFFFD; (*aktu&#xFFFD; (*aktu&#xFFFD; (*aktu&#xFFFD; (*aktu&#xFFFD; (*aktu&#xFFFD; (*aktu&#xFFFD; (*aktu&#xFFFD; (*aktu&#xFFFD; (*aktu&#xFFFD; (*aktu&#xFFFD; (*aktu&#xFFFD; (*aktu&#xFFFD; (*aktu&#xFFFD; (*aktu&#xFFFD; (*aktu&#xFFFD; (*aktu&#xFFFD; (*aktu&#xFFFD; (*aktu&#xFFFD; (*aktu&#xFFFD; (*aktu&#xFFFD; (*aktu&#xFFFD; (*aktu&#xFFFD; (*aktu&#xFFFD; (*aktu&#xFFFD; (*aktu&#xFFFD; (*aktu&#xFFFD; (*aktu&#xFFFD; (*aktu&#xFFFD; (*aktu&#xFFFD; (*aktu&#xFFFD; (*aktu&#xFFFD; (*aktu&#xFFFD; (*aktu&#xFFFD; (*aktu&#xFFFD; (*aktu&#xFFFD; (*aktu&#xFFFD; (*aktu&#xFFFD; (*aktu&#xFFFD; (*aktu&#xFFFD; (*aktu&#xFFFD; (*aktu&#xFFFD; (*aktu&#xFFFD; (*aktu&#xFFFD; (*aktu&#xFFFD; (*aktu&#xFFFD; (*aktu&#xFFFD; (*aktu&#xFFFD; (*aktu&#xFFFD; (*aktu&#xFFFD; (*aktu&#xFFFD; (*aktu&#xFFFD; (*aktu&#xFFFD; (*aktu&#xFFFD; (*aktu&#xFFFD; (*aktu&#xFFFD; (*aktu&#xFFFD; (*aktu&#xFFFD; (*aktu&#xFFFD; (*aktu&#xFFFD; (*aktu&#xFFFD; (*aktu&#xFFFD; (*aktu&#xFFFD; (*aktu&#xFFFD; (*aktu&#xFFFD; (*aktu&#xFFFD; (*aktu&#xFFFD; (*aktu&#xFFFD; (*aktu&#xFFFD; (*aktu&#xFFFD; (*aktu&#xFFFD; (*aktu&#xFFFD; (*aktu&#xFFFD; (*aktu&#xFFFD; (*aktu&#xFFFD; (*aktu&#xFFFD; (*aktu&#xFFFD; (*aktu&#xFFFD; (*aktu&#xFFFD; (*aktu&#xFFFD; (*aktu&#xFFFD; (*aktu&#xFFFD; (*aktu&#xFFFD; (*aktu&#xFFFD; (*aktu&#xFFFD; (*aktu&#xFFFD; (*aktu&#xFFFD; (*aktu&#xFFFD; (*aktu&#xFFFD; (*aktu&#xFFFD; (*aktu&#xFFFD; (*aktu&#xFFFD; (*aktu&#xFFFD; (*aktu&#xFFFD; (*aktu&#xFFFD; (*aktu&#xFFFD; (*aktu&#xFFFD; (*aktu&#xFFFD; (*aktu&#xFFFD; (*aktu&#xFFFD; (*aktu&#xFFFD; (*aktu&#xFFFD; (*aktu&#xFFFD; (*aktu&#xFFFD; (*aktu&#xFFFD; (*aktu&#xFFFD; (*aktu&#xFFFD; (*aktu&#xFFFD; (*aktu&#xFFFD; (*aktu&#xFFFD; (*aktu&#xFFFD; (*aktu&#xFFFD; (*aktu&#xFFFD; (*aktu&#xFFFD; (*aktu&#xFFFD; (*aktu&#xFFFD; (*aktu&#xFFFD; (*aktu&#xFFFD; (*aktu&#xFFFD; (*aktu&#xFFFD; (*aktu&#xFFFD; (*aktu&#xFFFD; (*aktu&#xFFFD; (*aktu&#xFFFD; (*aktu&#xFFFD; (*aktu&#xFFFD; (*aktu&#xFFFD; (*aktu&#xFFFD; (*aktu&#xFFFD; (*aktu&#xFFFD; (*aktu&#xFFFD; (*aktu&#xFFFD; (*aktu&#xFFFD; (*aktu&#xFFFD; (*aktu&#xFFFD; (*aktu&#xFFFD; (*aktu&#xFFFD; (*aktu&#xFFFD; (*aktu&#xFFFD; (*aktu&#xFFFD; (*aktu&#xFFFD; (*aktu&#xFFFD; (*aktu&#xFFFD; (*aktu&#xFFFD; (*aktu&#xFFFD; (*aktu&#xFFFD; (*aktu&#xFFFD; (*aktu&#xFFFD; (*aktu&#xFFFD; (*aktu&#xFFFD; (*aktu&#xFFFD; (*aktu&#xFFFD; (*aktu&#xFFFD; (*aktu&#xFFFD; (*aktu&#xFFFD; (*aktu&#xFFFD; (*aktu&#xFFFD; (*aktu&#xFFFD; (*aktu&#xFFFD; (*aktu&#xFFFD; (*aktu&#xFFFD; (*aktu&#xFFFD; (*aktu&#xFFFD; (*aktu&#xFFFD; (*aktu&#xFFFD; (*aktu&#xFFFD; (*aktu&#xFFFD; (*aktu&#xFFFD; (*aktu&#xFFFD; (*aktu&#xFFFD; (*aktu&#xFFFD; (*aktu&#xFFFD; (*aktu&#xFFFD; (*aktu&#xFFFD; (*aktu&#xFFFD; (*aktu&#xFFFD; (*aktu&#xFFFD; (*aktu&#xFFFD; (*aktu&#xFFFD; (*aktu&#xFFFD; (*aktu&#xFFFD; (*aktu&#xFFFD; (*aktu&#xFFFD; (*aktu&#xFFFD; (*aktu&#xFFFD; (*aktu&#xFFFD; (*aktu&#xFFFD; (*aktu&#xFFFD; (*aktu&#xFFFD; (*aktu&#xFFFD; (*aktu&#xFFFD; (*aktu&#xFFFD; (*aktu&#xFFFD; (*aktu&#xFFFD; (*aktu&#xFFFD; (*aktu&#xFFFD; (*aktu&#xFFFD; (*aktu&#xFFFD; (*aktu&#xFFFD; (*aktu&#xFFFD; (*aktu&#xFFFD; (*aktu&#xFFFD; (*aktu&#xFFFD; (*aktu&#xFFFD; (*aktu&#xFFFD; (*aktu&#xFFFD; (*aktu&#xFFFD; (*aktu&#xFFFD; (*aktu&#xFFFD; (*aktu&#xFFFD; (*aktu&#xFFFD; (*aktu&#xFFFD; (*aktu&#xFFFD; (*aktu&#xFFFD; (*aktu&#xFFFD; (*aktu&#xFFFD; (*aktu&#xFFFD; (*aktu&#xFFFD; (*aktu&#xFFFD; (*aktu&#xFFFD; (*aktu&#xFFFD; (*aktu&#xFFFD; (*aktu&#xFFFD; (*aktu&#xFFFD; (*aktu&#xFFFD; (*aktu&#xFFFD; (*aktu&#xFFFD; (*aktu&#xFFFD; (*aktu&#xFFFD; (*aktu&#xFFFD; (*aktu&#xFFFD; (*aktu&#xFFFD; (*aktu&#xFFFD; (*aktu&#xFFFD; (*aktu&#xFFFD; (*aktu&#xFFFD; (*aktu&#xFFFD; (*aktu&#xFFFD; (*aktu&#xFFFD; (*aktu&#xFFFD; (*aktu&#xFFFD; (*aktu&#xFFFD; (*aktu&#xFFFD; (*aktu&#xFFFD; (*aktu&#xFFFD; (*aktu&#xFFFD; (*aktu&#xFFFD; (*aktu&#xFFFD; (*aktu&#xFFFD; (*aktu&#xFFFD; (*aktu&#xFFFD; (*aktu&#xFFFD; (*aktu&#xFFFD; (*aktu&#xFFFD; (*aktu&#xFFFD; (*aktu&#xFFFD; (*aktu&#xFFFD; (*aktu&#xFFFD; (*aktu&#xFFFD; (*aktu&#xFFFD; (*aktu&#xFFFD; (*aktu&#xFFFD; (*aktu&#xFFFD; (*aktu&#xFFFD; (*aktu&#xFFFD; (*aktu&#xFFFD; (*aktu&#xFFFD; (*aktu&#xFFFD; (*aktu&#xFFFD; (*aktu&#xFFFD; (*aktu&#xFFFD; (*aktu&#xFFFD; (*aktu&#xFFFD; (*aktu&#xFFFD; (*aktu&#xFFFD; (*aktu&#xFFFD; (*aktu&#xFFFD; (*aktu&#xFFFD; (*aktu&#xFFFD; (*aktu&#xFFFD; (*aktu&#xFFFD; (*aktu&#xFFFD; (*aktu&#xFFFD; (*aktu&#xFFFD; (*aktu&#xFFFD; (*aktu&#xFFFD; (*aktu&#xFFFD; (*aktu&#xFFFD; (*aktu&#xFFFD; (*aktu&#xFFFD; (*aktu&#xFFFD; (*aktu&#xFFFD; (*aktu&#xFFFD; (*aktu&#xFFFD; (*aktu&#xFFFD; (*aktu&#xFFFD; (*aktu&#xFFFD; (*aktu&#xFFFD; (*aktu&#xFFFD; (*aktu&#xFFFD; (*aktu&#xFFFD; (*aktu&#xFFFD; (*aktu&#xFFFD; (*aktu&#xFFFD; (*aktu&#xFFFD; (*aktu&#xFFFD; (*aktu&#xFFFD; (*aktu&#xFFFD; (*aktu&#xFFFD; (*aktu&#xFFFD; (*aktu&#xFFFD; (*aktu&#xFFFD; (*aktu&#xFFFD; (*aktu&#xFFFD; (*aktu&#xFFFD; (*aktu&#xFFFD; (*aktu&#xFFFD; (*aktu&#xFFFD; (*aktu&#xFFFD; (*aktu&#xFFFD; (*aktu&#xFFFD; (*aktu&#xFFFD; (*aktu&#xFFFD; (*aktu&#xFFFD; (*aktu&#xFFFD; (*aktu&#xFFFD; (*aktu&#xFFFD; (*aktu&#xFFFD; (*aktu&#xFFFD; (*aktu&#xFFFD; (*aktu&#xFFFD; (*aktu&#xFFFD; (*aktu&#xFFFD; (*aktu&#xFFFD; (*aktu&#xFFFD; (*aktu&#xFFFD; (*aktu&#xFFFD; (*aktu&#xFFFD; (*aktu&#xFFFD; (*aktu&#xFFFD; (*aktu&#xFFFD; (*aktu&#xFFFD; (*aktu&#xFFFD; (*aktu&#xFFFD; (*aktu&#xFFFD; (*aktu&#xFFFD; (*aktu&#xFFFD; (*aktu&#xFFFD; (*aktu&#xFFFD; (*aktu&#xFFFD; (*aktu&#xFFFD; (*aktu&#xFFFD; (*aktu&#xFFFD; (*aktu&#xFFFD; (*aktu&#xFFFD; (*aktu&#xFFFD; (*aktu&#xFFFD; (*aktu&#xFFFD; (*aktu&#xFFFD; (*aktu&#xFFFD; (*aktu&#xFFFD; (*aktu&#xFFFD; (*aktu&#xFFFD; (*aktu&#xFFFD; (*aktu&#xFFFD; (*aktu&#xFFFD; (*aktu&#xFFFD; (*aktu&#xFFFD; (*aktu&#xFFFD; (*aktu&#xFFFD; (*aktu&#xFFFD; (*aktu&#xFFFD; (*aktu&#xFFFD; (*aktu&#xFFFD; (*aktu&#xFFFD; (*aktu&#xFFFD; (*aktu&#xFFFD; (*aktu&#xFFFD; (*aktu&#xFFFD; (*aktu&#xFFFD; (*aktu&#xFFFD; (*aktu&#xFFFD; (*aktu&#xFFFD; (*aktu&#xFFFD; (*aktu&#xFFFD; (*aktu&#xFFFD; (*aktu&#xFFFD; (*aktu&#xFFFD; (*aktu&#xFFFD; (*aktu&#xFFFD; (*aktu&#xFFFD; (*aktu&#xFFFD; (*aktu&#xFFFD; (*aktu&#xFFFD; (*aktu&#xFFFD; (*aktu&#xFFFD; (*aktu&#xFFFD; (*aktu&#xFFFD; (*aktu&#xFFFD; (*aktu&#xFFFD; (*aktu&#xFFFD; (*aktu&#xFFFD; (*aktu&#xFFFD; (*aktu&#xFFFD; (*aktu&#xFFFD; (*aktu&#xFFFD; (*aktu&#xFFFD; (*aktu&#xFFFD; (*aktu&#xFFFD; (*aktu&#xFFFD; (*aktu&#xFFFD; (*aktu&#xFFFD; (*aktu&#xFFFD; (*aktu&#xFFFD; (*aktu&#xFFFD; (*aktu&#xFFFD; (*aktu&#xFFFD; (*aktu&#xFFFD; (*aktu&#xFFFD; (*aktu&#xFFFD; (*aktu&#xFFFD; (*aktu&#xFFFD; (*aktu&#xFFFD; (*aktu&#xFFFD; (*aktu&#xFFFD; (*aktu&#xFFFD; (*aktu&#xFFFD; (*aktu&#xFFFD; (*aktu&#xFFFD; (*aktu&#xFFFD; (*aktu&#xFFFD; (*aktu&#xFFFD; (*aktu&#xFFFD; (*aktu&#xFFFD; (*aktu&#xFFFD; (*aktu&#xFFFD; (*aktu&#xFFFD; (*aktu&#xFFFD; (*aktu&#xFFFD; (*aktu&#xFFFD; (*aktu&#xFFFD; (*aktu&#xFFFD; (*aktu&#xFFFD; (*aktu&#xFFFD; (*aktu&#xFFFD; (*aktu&#xFFFD; (*aktu&#xFFFD; (*aktu&#xFFFD; (*aktu&#xFFFD; (*aktu&#xFFFD; (*aktu&#xFFFD; (*aktu&#xFFFD; (*aktu&#xFFFD; (*aktu&#xFFFD; (*aktu&#xFFFD; (*aktu&#xFFFD; (*aktu&#xFFFD; (*aktu&#xFFFD; (*aktu&#xFFFD; (*aktu&#xFFFD; (*aktu&#xFFFD; (*aktu&#xFFFD; (*aktu&#xFFFD; (*aktu&#xFFFD; (*aktu&#xFFFD; (*aktu&#xFFFD; (*aktu&#xFFFD; (*aktu&#xFFFD; (*aktu&#xFFFD; (*aktu&#xFFFD; (*aktu&#xFFFD; (*aktu&#xFFFD; (*aktu&#xFFFD; (*aktu&#xFFFD; (*aktu&#xFFFD; (*aktu&#xFFFD; (*aktu&#xFFFD; (*aktu&#xFFFD; (*aktu&#xFFFD; (*aktu&#xFFFD; (*aktu&#xFFFD; (*aktu&#xFFFD; (*aktu&#xFFFD; (*aktu&#xFFFD; (*aktu&#xFFFD; (*aktu&#xFFFD; (*aktu&#xFFFD; (*aktu&#xFFFD; (*aktu&#xFFFD; (*aktu&#xFFFD; (*aktu&#xFFFD; (*aktu&#xFFFD; (*aktu&#xFFFD; (*aktu&#xFFFD; (*aktu&#xFFFD; (*aktu&#xFFFD; (*aktu&#xFFFD; (*aktu&#xFFFD; (*aktu&#xFFFD; (*aktu&#xFFFD; (*aktu&#xFFFD; (*aktu&#xFFFD; (*aktu&#xFFFD; (*aktu&#xFFFD; (*aktu&#xFFFD; (*aktu&#xFFFD; (*aktu&#xFFFD; (*aktu&#xFFFD; (*aktu&#xFFFD; (*aktu&#xFFFD; (*aktu&#xFFFD; (*aktu&#xFFFD; (*aktu&#xFFFD; (*aktu&#xFFFD; (*aktu&#xFFFD; (*aktu&#xFFFD; (*aktu&#xFFFD; (*aktu&#xFFFD; (*aktu&#xFFFD; (*aktu&#xFFFD; (*aktu&#xFFFD; (*aktu&#xFFFD; (*aktu&#xFFFD; (*aktu&#xFFFD; (*aktu&#xFFFD; (*aktu&#xFFFD; (*aktu&#xFFFD; (*aktu&#xFFFD; (*aktu&#xFFFD; (*aktu&#xFFFD; (*aktu&#xFFFD; (*aktu&#xFFFD; (*aktu&#xFFFD; (*aktu&#xFFFD; (*aktu&#xFFFD; (*aktu&#xFFFD; (*aktu&#xFFFD; (*aktu&#xFFFD; (*aktu&#xFFFD; (*aktu&#xFFFD; (*aktu&#xFFFD; (*aktu&#xFFFD; (*aktu&#xFFFD; (*aktu&#xFFFD; (*aktu&#xFFFD; (*aktu&#xFFFD; (*aktu&#xFFFD; (*aktu&#xFFFD; (*aktu&#xFFFD; (*aktu&#xFFFD; (*aktu&#xFFFD; (*aktu&#xFFFD; (*aktu&#xFFFD; (*aktu&#xFFFD; (*aktu&#xFFFD; (*aktu&#xFFFD; (*aktu&#xFFFD; (*aktu&#xFFFD; (*aktu&#xFFFD; (*aktu&#xFFFD; (*aktu&#xFFFD; (*aktu&#xFFFD; (*aktu&#xFFFD; (*aktu&#xFFFD; (*aktu&#xFFFD; (*aktu&#xFFFD; (*aktu&#xFFFD; (*aktu&#xFFFD; (*aktu&#xFFFD; (*aktu&#xFFFD; (*aktu&#xFFFD; (*aktu&#xFFFD; (*aktu&#xFFFD; (*aktu&#xFFFD; (*aktu&#xFFFD; (*aktu&#xFFFD; (*aktu&#xFFFD; (*aktu&#xFFFD; (*aktu&#xFFFD; (*aktu&#xFFFD; (*aktu&#xFFFD; (*aktu&#xFFFD; (*aktu&#xFFFD; (*aktu&#xFFFD; (*aktu&#xFFFD; (*aktu&#xFFFD; (*aktu&#xFFFD; (*aktu&#xFFFD; (*aktu&#xFFFD; (*aktu&#xFFFD; (*aktu&#xFFFD; (*aktu&#xFFFD; (*aktu&#xFFFD; (*aktu&#xFFFD; (*aktu&#xFFFD; (*aktu&#xFFFD; (*aktu&#xFFFD; (*aktu&#xFFFD; (*aktu&#xFFFD; (*aktu&#xFFFD; (*aktu&#xFFFD; (*aktu&#xFFFD; (*aktu&#xFFFD; (*aktu&#xFFFD; (*aktu&#xFFFD; (*aktu&#xFFFD; (*aktu&#xFFFD; (*aktu&#xFFFD; (*aktu&#xFFFD; (*aktu&#xFFFD; (*aktu&#xFFFD; (*aktu&#xFFFD; (*aktu&#xFFFD; (*aktu&#xFFFD; (*aktu&#xFFFD; (*aktu&#xFFFD; (*aktu&#xFFFD; (*aktu&#xFFFD; (*aktu&#xFFFD; (*aktu&#xFFFD; (*aktu&#xFFFD; (*aktu&#xFFFD; (*aktu&#xFFFD; (*aktu&#xFFFD; (*aktu&#xFFFD; (*aktu&#xFFFD; (*aktu&#xFFFD; (*aktu&#xFFFD; (*aktu&#xFFFD; (*aktu&#xFFFD; (*aktu&#xFFFD; (*aktu&#xFFFD; (*aktu&#xFFFD; (*aktu&#xFFFD; (*aktu&#xFFFD; (*aktu&#xFFFD; (*aktu&#xFFFD; (*aktu&#xFFFD; (*aktu&#xFFFD; (*aktu&#xFFFD; (*aktu&#xFFFD; (*aktu&#xFFFD; (*aktu&#xFFFD; (*aktu&#xFFFD; (*aktu&#xFFFD; (*aktu&#xFFFD; (*aktu&#xFFFD; (*aktu&#xFFFD; (*aktu&#xFFFD; (*aktu&#xFFFD; (*aktu&#xFFFD; (*aktu&#xFFFD; (*aktu&#xFFFD; (*aktu&#xFFFD; (*aktu&#xFFFD; (*aktu&#xFFFD; (*aktu&#xFFFD; (*aktu&#xFFFD; (*aktu&#xFFFD; (*aktu&#xFFFD; (*aktu&#xFFFD; (*aktu&#xFFFD; (*aktu&#xFFFD; (*aktu&#xFFFD; (*aktu&#xFFFD; (*aktu&#xFFFD; (*aktu&#xFFFD; (*aktu&#xFFFD; (*aktu&#xFFFD; (*aktu&#xFFFD; (*aktu&#xFFFD; (*aktu&#xFFFD; (*aktu&#xFFFD; (*aktu&#xFFFD; (*aktu&#xFFFD; (*aktu&#xFFFD; (*aktu&#xFFFD; (*aktu&#xFFFD; (*aktu&#xFFFD; (*aktu&#xFFFD; (*aktu&#xFFFD; (*aktu&#xFFFD; (*aktu&#xFFFD; (*aktu&#xFFFD; (*aktu&#xFFFD; (*aktu&#xFFFD; (*aktu&#xFFFD; (*aktu&#xFFFD; (*aktu&#xFFFD; (*aktu&#xFFFD; (*aktu&#xFFFD; (*aktu&#xFFFD; (*aktu&#xFFFD; (*aktu&#xFFFD; (*aktu&#xFFFD; (*aktu&#xFFFD; (*aktu&#xFFFD; (*aktu&#xFFFD; (*aktu&#xFFFD; (*aktu&#xFFFD; (*aktu&#xFFFD; (*aktu&#xFFFD; (*aktu&#xFFFD; (*aktu&#xFFFD; (*aktu&#xFFFD; (*aktu&#xFFFD; (*aktu&#xFFFD; (*aktu&#xFFFD; (*aktu&#xFFFD; (*aktu&#xFFFD; (*aktu&#xFFFD; (*aktu&#xFFFD; (*aktu&#xFFFD; (*aktu&#xFFFD; (*aktu&#xFFFD; (*aktu&#xFFFD; (*aktu&#xFFFD; (*aktu&#xFFFD; (*aktu&#xFFFD; (*aktu&#xFFFD; (*aktu&#xFFFD; (*aktu&#xFFFD; (*aktu&#xFFFD; (*aktu&#xFFFD; (*aktu&#xFFFD; (*aktu&#xFFFD; (*aktu&#xFFFD; (*aktu&#xFFFD; (*aktu&#xFFFD; (*aktu&#xFFFD; (*aktu&#xFFFD; (*aktu&#xFFFD; (*aktu&#xFFFD; (*aktu&#xFFFD; (*aktu&#xFFFD; (*aktu&#xFFFD; (*aktu&#xFFFD; (*aktu&#xFFFD; (*aktu&#xFFFD; (*aktu&#xFFFD; (*aktu&#xFFFD; (*aktu&#xFFFD; (*aktu&#xFFFD; (*aktu&#xFFFD; (*aktu&#xFFFD; (*aktu&#xFFFD; (*aktu&#xFFFD; (*aktu&#xFFFD; (*aktu&#xFFFD; (*aktu&#xFFFD; (*aktu&#xFFFD; (*aktu&#xFFFD; (*aktu&#xFFFD; (*aktu&#xFFFD; (*aktu&#xFFFD; (*aktu&#xFFFD; (*aktu&#xFFFD; (*aktu&#xFFFD; (*aktu&#xFFFD; (*aktu&#xFFFD; (*aktu&#xFFFD; (*aktu&#xFFFD; (*aktu&#xFFFD; (*aktu&#xFFFD; (*aktu&#xFFFD; (*aktu&#xFFFD; (*aktu&#xFFFD; (*aktu&#xFFFD; (*aktu&#xFFFD; (*aktu&#xFFFD; (*aktu&#xFFFD; (*aktu&#xFFFD; (*aktu&#xFFFD; (*aktu&#xFFFD; (*aktu&#xFFFD; (*aktu&#xFFFD; (*aktu&#xFFFD; (*aktu&#xFFFD; (*aktu&#xFFFD; (*aktu&#xFFFD; (*aktu&#xFFFD; (*aktu&#xFFFD; (*aktu&#xFFFD; (*aktu&#xFFFD; (*aktu&#xFFFD; (*aktu&#xFFFD; (*aktu&#xFFFD; (*aktu&#xFFFD; (*aktu&#xFFFD; (*aktu&#xFFFD; (*aktu&#xFFFD; (*aktu&#xFFFD; (*aktu&#xFFFD; (*aktu&#xFFFD; (*aktu&#xFFFD; (*aktu&#xFFFD; (*aktu&#xFFFD; (*aktu&#xFFFD; (*aktu&#xFFFD; (*aktu&#xFFFD; (*aktu&#xFFFD; (*aktu&#xFFFD; (*aktu&#xFFFD; (*aktu&#xFFFD; (*aktu&#xFFFD; (*aktu&#xFFFD; (*aktu&#xFFFD; (*aktu&#xFFFD; (*aktu&#xFFFD; (*aktu&#xFFFD; (*aktu&#xFFFD; (*aktu&#xFFFD; (*aktu&#xFFFD; (*aktu&#xFFFD; (*aktu&#xFFFD; (*aktu&#xFFFD; (*aktu&#xFFFD; (*aktu&#xFFFD; (*aktu&#xFFFD; (*aktu&#xFFFD; (*aktu&#xFFFD; (*aktu&#xFFFD; (*aktu&#xFFFD; (*aktu&#xFFFD; (*aktu&#xFFFD; (*aktu&#xFFFD; (*aktu&#xFFFD; (*aktu&#xFFFD; (*aktu&#xFFFD; (*aktu&#xFFFD; (*aktu&#xFFFD; (*aktu&#xFFFD; (*aktu&#xFFFD; (*aktu&#xFFFD; (*aktu&#xFFFD; (*aktu&#xFFFD; (*aktu&#xFFFD; (*aktu&#xFFFD; (*aktu&#xFFFD; (*aktu&#xFFFD; (*aktu&#xFFFD; (*aktu&#xFFFD; (*aktu&#xFFFD; (*aktu&#xFFFD; (*aktu&#xFFFD; (*aktu&#xFFFD; (*aktu&#xFFFD; (*aktu&#xFFFD; (*aktu&#xFFFD; (*aktu&#xFFFD; (*aktu&#xFFFD; (*aktu&#xFFFD; (*aktu&#xFFFD; (*aktu&#xFFFD; (*aktu&#xFFFD; (*aktu&#xFFFD; (*aktu&#xFFFD; (*aktu&#xFFFD; (*aktu&#xFFFD; (*aktu&#xFFFD; (*aktu&#xFFFD; (*aktu&#xFFFD; (*aktu&#xFFFD; (*aktu&#xFFFD; (*aktu&#xFFFD; (*aktu&#xFFFD; (*aktu&#xFFFD; (*aktu&#xFFFD; (*aktu&#xFFFD; (*aktu&#xFFFD; (*aktu&#xFFFD; (*aktu&#xFFFD; (*aktu&#xFFFD; (*aktu&#xFFFD; (*aktu&#xFFFD; (*aktu&#xFFFD; (*aktu&#xFFFD; (*aktu&#xFFFD; (*aktu&#xFFFD; (*aktu&#xFFFD; (*aktu&#xFFFD; (*aktu&#xFFFD; (*aktu&#xFFFD; (*aktu&#xFFFD; (*aktu&#xFFFD; (*aktu&#xFFFD; (*aktu&#xFFFD; (*aktu&#xFFFD; (*aktu&#xFFFD; (*aktu&#xFFFD; (*aktu&#xFFFD; (*aktu&#xFFFD; (*aktu&#xFFFD; (*aktu&#xFFFD; (*aktu&#xFFFD; (*aktu&#xFFFD; (*aktu&#xFFFD; (*aktu&#xFFFD; (*aktu&#xFFFD; (*aktu&#xFFFD; (*aktu&#xFFFD; (*aktu&#xFFFD; (*aktu&#xFFFD; (*aktu&#xFFFD; (*aktu&#xFFFD; (*aktu&#xFFFD; (*aktu&#xFFFD; (*aktu&#xFFFD; (*aktu&#xFFFD; (*aktu&#xFFFD; (*aktu&#xFFFD; (*aktu&#xFFFD; (*aktu&#xFFFD; (*aktu&#xFFFD; (*aktu&#xFFFD; (*aktu&#xFFFD; (*aktu&#xFFFD; (*aktu&#xFFFD; (*aktu&#xFFFD; (*aktu&#xFFFD; (*aktu&#xFFFD; (*aktu&#xFFFD; (*aktu&#xFFFD; (*aktu&#xFFFD; (*aktu&#xFFFD; (*aktu&#xFFFD; (*aktu&#xFFFD; (*aktu&#xFFFD; (*aktu&#xFFFD; (*aktu&#xFFFD; (*aktu&#xFFFD; (*aktu&#xFFFD; (*aktu&#xFFFD; (*aktu&#xFFFD; (*aktu&#xFFFD; (*aktu&#xFFFD; (*aktu&#xFFFD; (*aktu&#xFFFD; (*aktu&#xFFFD; (*aktu&#xFFFD; (*aktu&#xFFFD; (*aktu&#xFFFD; (*aktu&#xFFFD; (*aktu&#xFFFD; (*aktu&#xFFFD; (*aktu&#xFFFD; (*aktu&#xFFFD; (*aktu&#xFFFD; (*aktu&#xFFFD; (*aktu&#xFFFD; (*aktu&#xFFFD; (*aktu&#xFFFD; (*aktu&#xFFFD; (*aktu&#xFFFD; (*aktu&#xFFFD; (*aktu&#xFFFD; (*aktu&#xFFFD; (*aktu&#xFFFD; (*aktu&#xFFFD; (*aktu&#xFFFD; (*aktu&#xFFFD; (*aktu&#xFFFD; (*aktu&#xFFFD; (*aktu&#xFFFD; (*aktu&#xFFFD; (*aktu&#xFFFD; (*aktu&#xFFFD; (*aktu&#xFFFD; (*aktu&#xFFFD; (*aktu&#xFFFD; (*aktu&#xFFFD; (*aktu&#xFFFD; (*aktu&#xFFFD; (*aktu&#xFFFD; (*aktu&#xFFFD; (*aktu&#xFFFD; (*aktu&#xFFFD; (*aktu&#xFFFD; (*aktu&#xFFFD; (*aktu&#xFFFD; (*aktu&#xFFFD; (*aktu&#xFFFD; (*aktu&#xFFFD; (*aktu&#xFFFD; (*aktu&#xFFFD; (*aktu&#xFFFD; (*aktu&#xFFFD; (*aktu&#xFFFD; (*aktu&#xFFFD; (*aktu&#xFFFD; (*aktu&#xFFFD; (*aktu&#xFFFD; (*aktu&#xFFFD; (*aktu&#xFFFD; (*aktu&#xFFFD; (*aktu&#xFFFD; (*aktu&#xFFFD; (*aktu&#xFFFD; (*aktu&#xFFFD; (*aktu&#xFFFD; (*aktu&#xFFFD; (*aktu&#xFFFD; (*aktu&#xFFFD; (*aktu&#xFFFD; (*aktu&#xFFFD; (*aktu&#xFFFD; (*aktu&#xFFFD; (*aktu&#xFFFD; (*aktu&#xFFFD; (*aktu&#xFFFD; (*aktu&#xFFFD; (*aktu&#xFFFD; (*aktu&#xFFFD; (*aktu&#xFFFD; (*aktu&#xFFFD; (*aktu&#xFFFD; (*aktu&#xFFFD; (*aktu&#xFFFD; (*aktu&#xFFFD; (*aktu&#xFFFD; (*aktu&#xFFFD; (*aktu&#xFFFD; (*aktu&#xFFFD; (*aktu&#xFFFD; (*aktu&#xFFFD; (*aktu&#xFFFD; (*aktu&#xFFFD; (*aktu&#xFFFD; (*aktu&#xFFFD; (*aktu&#xFFFD; (*aktu&#xFFFD; (*aktu&#xFFFD; (*aktu&#xFFFD; (*aktu&#xFFFD; (*aktu&#xFFFD; (*aktu&#xFFFD; (*aktu&#xFFFD; (*aktu&#xFFFD; (*aktu&#xFFFD; (*aktu&#xFFFD; (*aktu&#xFFFD; (*aktu&#xFFFD; (*aktu&#xFFFD; (*aktu&#xFFFD; (*aktu&#xFFFD; (*aktu&#xFFFD; (*aktu&#xFFFD; (*aktu&#xFFFD; (*aktu&#xFFFD; (*aktu&#xFFFD; (*aktu&#xFFFD; (*aktu&#xFFFD; (*aktu&#xFFFD; (*aktu&#xFFFD; (*aktu&#xFFFD; (*aktu&#xFFFD; (*aktu&#xFFFD; (*aktu&#xFFFD; (*aktu&#xFFFD; (*aktu&#xFFFD; (*aktu&#xFFFD; (*aktu&#xFFFD; (*aktu&#xFFFD; (*aktu&#xFFFD; (*aktu&#xFFFD; (*aktu&#xFFFD; (*aktu&#xFFFD; (*aktu&#xFFFD; (*aktu&#xFFFD; (*aktu&#xFFFD; (*aktu&#xFFFD; (*aktu&#xFFFD; (*aktu&#xFFFD; (*aktu&#xFFFD; (*aktu&#xFFFD; (*aktu&#xFFFD; (*aktu&#xFFFD; (*aktu&#xFFFD; (*aktu&#xFFFD; (*aktu&#xFFFD; (*aktu&#xFFFD; (*aktu&#xFFFD; (*aktu&#xFFFD; (*aktu&#xFFFD; (*aktu&#xFFFD; (*aktu&#xFFFD; (*aktu&#xFFFD; (*aktu&#xFFFD; (*aktu&#xFFFD; (*aktu&#xFFFD; (*aktu&#xFFFD; (*aktu&#xFFFD; (*aktu&#xFFFD; (*aktu&#xFFFD; (*aktu&#xFFFD; (*aktu&#xFFFD; (*aktu&#xFFFD; (*aktu&#xFFFD; (*aktu&#xFFFD; (*aktu&#xFFFD; (*aktu&#xFFFD; (*aktu&#xFFFD; (*aktu&#xFFFD; (*aktu&#xFFFD; (*aktu&#xFFFD; (*aktu&#xFFFD; (*aktu&#xFFFD; (*aktu&#xFFFD; (*aktu&#xFFFD; (*aktu&#xFFFD; (*aktu&#xFFFD; (*aktu&#xFFFD; (*aktu&#xFFFD; (*aktu&#xFFFD; (*aktu&#xFFFD; (*aktu&#xFFFD; (*aktu&#xFFFD; (*aktu&#xFFFD; (*aktu&#xFFFD; (*aktu&#xFFFD; (*aktu&#xFFFD; (*aktu&#xFFFD; (*aktu&#xFFFD; (*aktu&#xFFFD; (*aktu&#xFFFD; (*aktu&#xFFFD; (*aktu&#xFFFD; (*aktu&#xFFFD; (*aktu&#xFFFD; (*aktu&#xFFFD; (*aktu&#xFFFD; (*aktu&#xFFFD; (*aktu&#xFFFD; (*aktu&#xFFFD; (*aktu&#xFFFD; (*aktu&#xFFFD; (*aktu&#xFFFD; (*aktu&#xFFFD; (*aktu&#xFFFD; (*aktu&#xFFFD; (*aktu&#xFFFD; (*aktu&#xFFFD; (*aktu&#xFFFD; (*aktu&#xFFFD; (*aktu&#xFFFD; (*aktu&#xFFFD; (*aktu&#xFFFD; (*aktu&#xFFFD; (*aktu&#xFFFD; (*aktu&#xFFFD; (*aktu&#xFFFD; (*aktu&#xFFFD; (*aktu&#xFFFD; (*aktu&#xFFFD; (*aktu&#xFFFD; (*aktu&#xFFFD; (*aktu&#xFFFD; (*aktu&#xFFFD; (*aktu&#xFFFD; (*aktu&#xFFFD; (*aktu&#xFFFD; (*aktu&#xFFFD; (*aktu&#xFFFD; (*aktu&#xFFFD; (*aktu&#xFFFD; (*aktu&#xFFFD; (*aktu&#xFFFD; (*aktu&#xFFFD; (*aktu&#xFFFD; (*aktu&#xFFFD; (*aktu&#xFFFD; (*aktu&#xFFFD; (*aktu&#xFFFD; (*aktu&#xFFFD; (*aktu&#xFFFD; (*aktu&#xFFFD; (*aktu&#xFFFD; (*aktu&#xFFFD; (*aktu&#xFFFD; (*aktu&#xFFFD; (*aktu&#xFFFD; (*aktu&#xFFFD; (*aktu&#xFFFD; (*aktu&#xFFFD; (*aktu&#xFFFD; (*aktu&#xFFFD; (*aktu&#xFFFD; (*aktu&#xFFFD; (*aktu&#xFFFD; (*aktu&#xFFFD; (*aktu&#xFFFD; (*aktu&#xFFFD; (*aktu&#xFFFD; (*aktu&#xFFFD; (*aktu&#xFFFD; (*aktu&#xFFFD; (*aktu&#xFFFD; (*aktu&#xFFFD; (*aktu&#xFFFD; (*aktu&#xFFFD; (*aktu&#xFFFD; (*aktu&#xFFFD; (*aktu&#xFFFD; (*aktu&#xFFFD; (*aktu&#xFFFD; (*aktu&#xFFFD; (*aktu&#xFFFD; (*aktu&#xFFFD; (*aktu&#xFFFD; (*aktu&#xFFFD; (*aktu&#xFFFD; (*aktu&#xFFFD; (*aktu&#xFFFD; (*aktu&#xFFFD; (*aktu&#xFFFD; (*aktu&#xFFFD; (*aktu&#xFFFD; (*aktu&#xFFFD; (*aktu&#xFFFD; (*aktu&#xFFFD; (*aktu&#xFFFD; (*aktu&#xFFFD; (*aktu&#xFFFD; (*aktu&#xFFFD; (*aktu&#xFFFD; (*aktu&#xFFFD; (*aktu&#xFFFD; (*aktu&#xFFFD; (*aktu&#xFFFD; (*aktu&#xFFFD; (*aktu&#xFFFD; (*aktu&#xFFFD; (*aktu&#xFFFD; (*aktu&#xFFFD; (*aktu&#xFFFD; (*aktu&#xFFFD; (*aktu&#xFFFD; (*aktu&#xFFFD; (*aktu&#xFFFD; (*aktu&#xFFFD; (*aktu&#xFFFD; (*aktu&#xFFFD; (*aktu&#xFFFD; (*aktu&#xFFFD; (*aktu&#xFFFD; (*aktu&#xFFFD; (*aktu&#xFFFD; (*aktu&#xFFFD; (*aktu&#xFFFD; (*aktu&#xFFFD; (*aktu&#xFFFD; (*aktu&#xFFFD; (*aktu&#xFFFD; (*aktu&#xFFFD; (*aktu&#xFFFD; (*aktu&#xFFFD; (*aktu&#xFFFD; (*aktu&#xFFFD; (*aktu&#xFFFD; (*aktu&#xFFFD; (*aktu&#xFFFD; (*aktu&#xFFFD; (*aktu&#xFFFD; (*aktu&#xFFFD; (*aktu&#xFFFD; (*aktu&#xFFFD; (*aktu&#xFFFD; (*aktu&#xFFFD; (*aktu&#xFFFD; (*aktu&#xFFFD; (*aktu&#xFFFD; (*aktu&#xFFFD; (*aktu&#xFFFD; (*aktu&#xFFFD; (*aktu&#xFFFD; (*aktu&#xFFFD; (*aktu&#xFFFD; (*aktu&#xFFFD; (*aktu&#xFFFD; (*aktu&#xFFFD; (*aktu&#xFFFD; (*aktu&#xFFFD; (*aktu&#xFFFD; (*aktu&#xFFFD; (*aktu&#xFFFD; (*aktu&#xFFFD; (*aktu&#xFFFD; (*aktu&#xFFFD; (*aktu&#xFFFD; (*aktu&#xFFFD; (*aktu&#xFFFD; (*aktu&#xFFFD; (*aktu&#xFFFD; (*aktu&#xFFFD; (*aktu&#xFFFD; (*aktu&#xFFFD; (*aktu&#xFFFD; (*aktu&#xFFFD; (*aktu&#xFFFD; (*aktu&#xFFFD; (*aktu&#xFFFD; (*aktu&#xFFFD; (*aktu&#xFFFD; (*aktu&#xFFFD; (*aktu&#xFFFD; (*aktu&#xFFFD; (*aktu&#xFFFD; (*aktu&#xFFFD; (*aktu&#xFFFD; (*aktu&#xFFFD; (*aktu&#xFFFD; (*aktu&#xFFFD; (*aktu&#xFFFD; (*aktu&#xFFFD; (*aktu&#xFFFD; (*aktu&#xFFFD; (*aktu&#xFFFD; (*aktu&#xFFFD; (*aktu&#xFFFD; (*aktu&#xFFFD; (*aktu&#xFFFD; (*aktu&#xFFFD; (*aktu&#xFFFD; (*aktu&#xFFFD; (*aktu&#xFFFD; (*aktu&#xFFFD; (*aktu&#xFFFD; (*aktu&#xFFFD; (*aktu&#xFFFD; (*aktu&#xFFFD; (*aktu&#xFFFD; (*aktu&#xFFFD; (*aktu&#xFFFD; (*aktu&#xFFFD; (*aktu&#xFFFD; (*aktu&#xFFFD; (*aktu&#xFFFD; (*aktu&#xFFFD; (*aktu&#xFFFD; (*aktu&#xFFFD; (*aktu&#xFFFD; (*aktu&#xFFFD; (*aktu&#xFFFD; (*aktu&#xFFFD; (*aktu&#xFFFD; (*aktu&#xFFFD; (*aktu&#xFFFD; (*aktu&#xFFFD; (*aktu&#xFFFD; (*aktu&#xFFFD; (*aktu&#xFFFD; (*aktu&#xFFFD; (*aktu&#xFFFD; (*aktu&#xFFFD; (*aktu&#xFFFD; (*aktu&#xFFFD; (*aktu&#xFFFD; (*aktu&#xFFFD; (*aktu&#xFFFD; (*aktu&#xFFFD; (*aktu&#xFFFD; (*aktu&#xFFFD; (*aktu&#xFFFD; (*aktu&#xFFFD; (*aktu&#xFFFD; (*aktu&#xFFFD; (*aktu&#xFFFD; (*aktu&#xFFFD; (*aktu&#xFFFD; (*aktu&#xFFFD; (*aktu&#xFFFD; (*aktu&#xFFFD; (*aktu&#xFFFD; (*aktu&#xFFFD; (*aktu&#xFFFD; (*aktu&#xFFFD; (*aktu&#xFFFD; (*aktu&#xFFFD; (*aktu&#xFFFD; (*aktu&#xFFFD; (*aktu&#xFFFD; (*aktu&#xFFFD; (*aktu&#xFFFD; (*aktu&#xFFFD; (*aktu&#xFFFD; (*aktu&#xFFFD; (*aktu&#xFFFD; (*aktu&#xFFFD; (*aktu&#xFFFD; (*aktu&#xFFFD; (*aktu&#xFFFD; (*aktu&#xFFFD; (*aktu&#xFFFD; (*aktu&#xFFFD; (*aktu&#xFFFD; (*aktu&#xFFFD; (*aktu&#xFFFD; (*aktu&#xFFFD; (*aktu&#xFFFD; (*aktu&#xFFFD; (*aktu&#xFFFD; (*aktu&#xFFFD; (*aktu&#xFFFD; (*aktu&#xFFFD; (*aktu&#xFFFD; (*aktu&#xFFFD; (*aktu&#xFFFD; (*aktu&#xFFFD; (*aktu&#xFFFD; (*aktu&#xFFFD; (*aktu&#xFFFD; (*aktu&#xFFFD; (*aktu&#xFFFD; (*aktu&#xFFFD; (*aktu&#xFFFD; (*aktu&#xFFFD; (*aktu&#xFFFD; (*aktu&#xFFFD; (*aktu&#xFFFD; (*aktu&#xFFFD; (*aktu&#xFFFD; (*aktu&#xFFFD; (*aktu&#xFFFD; (*aktu&#xFFFD; (*aktu&#xFFFD; (*aktu&#xFFFD; (*aktu&#xFFFD; (*aktu&#xFFFD; (*aktu&#xFFFD; (*aktu&#xFFFD; (*aktu&#xFFFD; (*aktu&#xFFFD; (*aktu&#xFFFD; (*aktu&#xFFFD; (*aktu&#xFFFD; (*aktu&#xFFFD; (*aktu&#xFFFD; (*aktu&#xFFFD; (*aktu&#xFFFD; (*aktu&#xFFFD; (*aktu&#xFFFD; (*aktu&#xFFFD; (*aktu&#xFFFD; (*aktu&#xFFFD; (*aktu&#xFFFD; (*aktu&#xFFFD; (*aktu&#xFFFD; (*aktu&#xFFFD; (*aktu&#xFFFD; (*aktu&#xFFFD; (*aktu&#xFFFD; (*aktu&#xFFFD; (*aktu&#xFFFD; (*aktu&#xFFFD; (*aktu&#xFFFD; (*aktu&#xFFFD; (*aktu&#xFFFD; (*aktu&#xFFFD; (*aktu&#xFFFD; (*aktu&#xFFFD; (*aktu&#xFFFD; (*aktu&#xFFFD; (*aktu&#xFFFD; (*aktu&#xFFFD; (*aktu&#xFFFD; (*aktu&#xFFFD; (*aktu&#xFFFD; (*aktu&#xFFFD; (*aktu&#xFFFD; (*aktu&#xFFFD; (*aktu&#xFFFD; (*aktu&#xFFFD; (*aktu&#xFFFD; (*aktu&#xFFFD; (*aktu&#xFFFD; (*aktu&#xFFFD; (*aktu&#xFFFD; (*aktu&#xFFFD; (*aktu&#xFFFD; (*aktu&#xFFFD; (*aktu&#xFFFD; (*aktu&#xFFFD; (*aktu&#xFFFD; (*aktu&#xFFFD; (*aktu&#xFFFD; (*aktu&#xFFFD; (*aktu&#xFFFD; (*aktu&#xFFFD; (*aktu&#xFFFD; (*aktu&#xFFFD; (*aktu&#xFFFD; (*aktu&#xFFFD; (*aktu&#xFFFD; (*aktu&#xFFFD; (*aktu&#xFFFD; (*aktu&#xFFFD; (*aktu&#xFFFD; (*aktu&#xFFFD; (*aktu&#xFFFD; (*aktu&#xFFFD; (*aktu&#xFFFD; (*aktu&#xFFFD; (*aktu&#xFFFD; (*aktu&#xFFFD; (*aktu&#xFFFD; (*aktu&#xFFFD; (*aktu&#xFFFD; (*aktu&#xFFFD; (*aktu&#xFFFD; (*aktu&#xFFFD; (*aktu&#xFFFD; (*aktu&#xFFFD; (*aktu&#xFFFD; (*aktu&#xFFFD; (*aktu&#xFFFD; (*aktu&#xFFFD; (*aktu&#xFFFD; (*aktu&#xFFFD; (*aktu&#xFFFD; (*aktu&#xFFFD; (*aktu&#xFFFD; (*aktu&#xFFFD; (*aktu&#xFFFD; (*aktu&#xFFFD; (*aktu&#xFFFD; (*aktu&#xFFFD; (*aktu&#xFFFD; (*aktu&#xFFFD; (*aktu&#xFFFD; (*aktu&#xFFFD; (*aktu&#xFFFD; (*aktu&#xFFFD; (*aktu&#xFFFD; (*aktu&#xFFFD; (*aktu&#xFFFD; (*aktu&#xFFFD; (*aktu&#xFFFD; (*aktu&#xFFFD; (*aktu&#xFFFD; (*aktu&#xFFFD; (*aktu&#xFFFD; (*aktu&#xFFFD; (*aktu&#xFFFD; (*aktu&#xFFFD; (*aktu&#xFFFD; (*aktu&#xFFFD; (*aktu&#xFFFD; (*aktu&#xFFFD; (*aktu&#xFFFD; (*aktu&#xFFFD; (*aktu&#xFFFD; (*aktu&#xFFFD; (*aktu&#xFFFD; (*aktu&#xFFFD; (*aktu&#xFFFD; (*aktu&#xFFFD; (*aktu&#xFFFD; (*aktu&#xFFFD; (*aktu&#xFFFD; (*aktu&#xFFFD; (*aktu&#xFFFD; (*aktu&#xFFFD; (*aktu&#xFFFD; (*aktu&#xFFFD; (*aktu&#xFFFD; (*aktu&#xFFFD; (*aktu&#xFFFD; (*aktu&#xFFFD; (*aktu&#xFFFD; (*aktu&#xFFFD; (*aktu&#xFFFD; (*aktu&#xFFFD; (*aktu&#xFFFD; (*aktu&#xFFFD; (*aktu&#xFFFD; (*aktu&#xFFFD; (*aktu&#xFFFD; (*aktu&#xFFFD; (*aktu&#xFFFD; (*aktu&#xFFFD; (*aktu&#xFFFD; (*aktu&#xFFFD; (*aktu&#xFFFD; (*aktu&#xFFFD; (*aktu&#xFFFD; (*aktu&#xFFFD; (*aktu&#xFFFD; (*aktu&#xFFFD; (*aktu&#xFFFD; (*aktu&#xFFFD; (*aktu&#xFFFD; (*aktu&#xFFFD; (*aktu&#xFFFD; (*aktu&#xFFFD; (*aktu&#xFFFD; (*aktu&#xFFFD; (*aktu&#xFFFD; (*aktu&#xFFFD; (*aktu&#xFFFD; (*aktu&#xFFFD; (*aktu&#xFFFD; (*aktu&#xFFFD; (*aktu&#xFFFD; (*aktu&#xFFFD; (*aktu&#xFFFD; (*aktu&#xFFFD; (*aktu&#xFFFD; (*aktu&#xFFFD; (*aktu&#xFFFD; (*aktu&#xFFFD; (*aktu&#xFFFD; (*aktu&#xFFFD; (*aktu&#xFFFD; (*aktu&#xFFFD; (*aktu&#xFFFD; (*aktu&#xFFFD; (*aktu&#xFFFD; (*aktu&#xFFFD; (*aktu&#xFFFD; (*aktu&#xFFFD; (*aktu&#xFFFD; (*aktu&#xFFFD; (*aktu&#xFFFD; (*aktu&#xFFFD; (*aktu&#xFFFD; (*aktu&#xFFFD; (*aktu&#xFFFD; (*aktu&#xFFFD; (*aktu&#xFFFD; (*aktu&#xFFFD; (*aktu&#xFFFD; (*aktu&#xFFFD; (*aktu&#xFFFD; (*aktu&#xFFFD; (*aktu&#xFFFD; (*aktu&#xFFFD; (*aktu&#xFFFD; (*aktu&#xFFFD; (*aktu&#xFFFD; (*aktu&#xFFFD; (*aktu&#xFFFD; (*aktu&#xFFFD; (*aktu&#xFFFD; (*aktu&#xFFFD; (*aktu&#xFFFD; (*aktu&#xFFFD; (*aktu&#xFFFD; (*aktu&#xFFFD; (*aktu&#xFFFD; (*aktu&#xFFFD; (*aktu&#xFFFD; (*aktu&#xFFFD; (*aktu&#xFFFD; (*aktu&#xFFFD; (*aktu&#xFFFD; (*aktu&#xFFFD; (*aktu&#xFFFD; (*aktu&#xFFFD; (*aktu&#xFFFD; (*aktu&#xFFFD; (*aktu&#xFFFD; (*aktu&#xFFFD; (*aktu&#xFFFD; (*aktu&#xFFFD; (*aktu&#xFFFD; (*aktu&#xFFFD; (*aktu&#xFFFD; (*aktu&#xFFFD; (*aktu&#xFFFD; (*aktu&#xFFFD; (*aktu&#xFFFD; (*aktu&#xFFFD; (*aktu&#xFFFD; (*aktu&#xFFFD; (*aktu&#xFFFD; (*aktu&#xFFFD; (*aktu&#xFFFD; (*aktu&#xFFFD; (*aktu&#xFFFD; (*aktu&#xFFFD; (*aktu&#xFFFD; (*aktu&#xFFFD; (*aktu&#xFFFD; (*aktu&#xFFFD; (*aktu&#xFFFD; (*aktu&#xFFFD; (*aktu&#xFFFD; (*aktu&#xFFFD; (*aktu&#xFFFD; (*aktu&#xFFFD; (*aktu&#xFFFD; (*aktu&#xFFFD; (*aktu&#xFFFD; (*aktu&#xFFFD; (*aktu&#xFFFD; (*aktu&#xFFFD; (*aktu&#xFFFD; (*aktu&#xFFFD; (*aktu&#xFFFD; (*aktu&#xFFFD; (*aktu&#xFFFD; (*aktu&#xFFFD; (*aktu&#xFFFD; (*aktu&#xFFFD; (*aktu&#xFFFD; (*aktu&#xFFFD; (*aktu&#xFFFD; (*aktu&#xFFFD; (*aktu&#xFFFD; (*aktu&#xFFFD; (*aktu&#xFFFD; (*aktu&#xFFFD; (*aktu&#xFFFD; (*aktu&#xFFFD; (*aktu&#xFFFD; (*aktu&#xFFFD; (*aktu&#xFFFD; (*aktu&#xFFFD; (*aktu&#xFFFD; (*aktu&#xFFFD; (*aktu&#xFFFD; (*aktu&#xFFFD; (*aktu&#xFFFD; (*aktu&#xFFFD; (*aktu&#xFFFD; (*aktu&#xFFFD; (*aktu&#xFFFD; (*aktu&#xFFFD; (*aktu&#xFFFD; (*aktu&#xFFFD; (*aktu&#xFFFD; (*aktu&#xFFFD; (*aktu&#xFFFD; (*aktu&#xFFFD; (*aktu&#xFFFD; (*aktu&#xFFFD; (*aktu&#xFFFD; (*aktu&#xFFFD; (*aktu&#xFFFD; (*aktu&#xFFFD; (*aktu&#xFFFD; (*aktu&#xFFFD; (*aktu&#xFFFD; (*aktu&#xFFFD; (*aktu&#xFFFD; (*aktu&#xFFFD; (*aktu&#xFFFD; (*aktu&#xFFFD; (*aktu&#xFFFD; (*aktu&#xFFFD; (*aktu&#xFFFD; (*aktu&#xFFFD; (*aktu&#xFFFD; (*aktu&#xFFFD; (*aktu&#xFFFD; (*aktu&#xFFFD; (*aktu&#xFFFD; (*aktu&#xFFFD; (*aktu&#xFFFD; (*aktu&#xFFFD; (*aktu&#xFFFD; (*aktu&#xFFFD; (*aktu&#xFFFD; (*aktu&#xFFFD; (*aktu&#xFFFD; (*aktu&#xFFFD; (*aktu&#xFFFD; (*aktu&#xFFFD; (*aktu&#xFFFD; (*aktu&#xFFFD; (*aktu&#xFFFD; (*aktu&#xFFFD; (*aktu&#xFFFD; (*aktu&#xFFFD; (*aktu&#xFFFD; (*aktu&#xFFFD; (*aktu&#xFFFD; (*aktu&#xFFFD; (*aktu&#xFFFD; (*aktu&#xFFFD; (*aktu&#xFFFD; (*aktu&#xFFFD; (*aktu&#xFFFD; (*aktu&#xFFFD; (*aktu&#xFFFD; (*aktu&#xFFFD; (*aktu&#xFFFD; (*aktu&#xFFFD; (*aktu&#xFFFD; (*aktu&#xFFFD; (*aktu&#xFFFD; (*aktu&#xFFFD; (*aktu&#xFFFD; (*aktu&#xFFFD; (*aktu&#xFFFD; (*aktu&#xFFFD; (*aktu&#xFFFD; (*aktu&#xFFFD; (*aktu&#xFFFD; (*aktu&#xFFFD; (*aktu&#xFFFD; (*aktu&#xFFFD; (*aktu&#xFFFD; (*aktu&#xFFFD; (*aktu&#xFFFD; (*aktu&#xFFFD; (*aktu&#xFFFD; (*aktu&#xFFFD; (*aktu&#xFFFD; (*aktu&#xFFFD; (*aktu&#xFFFD; (*aktu&#xFFFD; (*aktu&#xFFFD; (*aktu&#xFFFD; (*aktu&#xFFFD; (*aktu&#xFFFD; (*aktu&#xFFFD; (*aktu&#xFFFD; (*aktu&#xFFFD; (*aktu&#xFFFD; (*aktu&#xFFFD; (*aktu&#xFFFD; (*aktu&#xFFFD; (*aktu&#xFFFD; (*aktu&#xFFFD; (*aktu&#xFFFD; (*aktu&#xFFFD; (*aktu&#xFFFD; (*aktu&#xFFFD; (*aktu&#xFFFD; (*aktu&#xFFFD; (*aktu&#xFFFD; (*aktu&#xFFFD; (*aktu&#xFFFD; (*aktu&#xFFFD; (*aktu&#xFFFD; (*aktu&#xFFFD; (*aktu&#xFFFD; (*aktu&#xFFFD; (*aktu&#xFFFD; (*aktu&#xFFFD; (*aktu&#xFFFD; (*aktu&#xFFFD; (*aktu&#xFFFD; (*aktu&#xFFFD; (*aktu&#xFFFD; (*aktu&#xFFFD; (*aktu&#xFFFD; (*aktu&#xFFFD; (*aktu&#xFFFD; (*aktu&#xFFFD; (*aktu&#xFFFD; (*aktu&#xFFFD; (*aktu&#xFFFD; (*aktu&#xFFFD; (*aktu&#xFFFD; (*aktu&#xFFFD; (*aktu&#xFFFD; (*aktu&#xFFFD; (*aktu&#xFFFD; (*aktu&#xFFFD; (*aktu&#xFFFD; (*aktu&#xFFFD; (*aktu&#xFFFD; (*aktu&#xFFFD; (*aktu&#xFFFD; (*aktu&#xFFFD; (*aktu&#xFFFD; (*aktu&#xFFFD; (*aktu&#xFFFD; (*aktu&#xFFFD; (*aktu&#xFFFD; (*aktu&#xFFFD; (*aktu&#xFFFD; (*aktu&#xFFFD; (*aktu&#xFFFD; (*aktu&#xFFFD; (*aktu&#xFFFD; (*aktu&#xFFFD; (*aktu&#xFFFD; (*aktu&#xFFFD; (*aktu&#xFFFD; (*aktu&#xFFFD; (*aktu&#xFFFD; (*aktu&#xFFFD; (*aktu&#xFFFD; (*aktu&#xFFFD; (*aktu&#xFFFD; (*aktu&#xFFFD; (*aktu&#xFFFD; (*aktu&#xFFFD; (*aktu&#xFFFD; (*aktu&#xFFFD; (*aktu&#xFFFD; (*aktu&#xFFFD; (*aktu&#xFFFD; (*aktu&#xFFFD; (*aktu&#xFFFD; (*aktu&#xFFFD; (*aktu&#xFFFD; (*aktu&#xFFFD; (*aktu&#xFFFD; (*aktu&#xFFFD; (*aktu&#xFFFD; (*aktu&#xFFFD; (*aktu&#xFFFD; (*aktu&#xFFFD; (*aktu&#xFFFD; (*aktu&#xFFFD; (*aktu&#xFFFD; (*aktu&#xFFFD; (*aktu&#xFFFD; (*aktu&#xFFFD; (*aktu&#xFFFD; (*aktu&#xFFFD; (*aktu&#xFFFD; (*aktu&#xFFFD; (*aktu&#xFFFD; (*aktu&#xFFFD; (*aktu&#xFFFD; (*aktu&#xFFFD; (*aktu&#xFFFD; (*aktu&#xFFFD; (*aktu&#xFFFD; (*aktu&#xFFFD; (*aktu&#xFFFD; (*aktu&#xFFFD; (*aktu&#xFFFD; (*aktu&#xFFFD; (*aktu&#xFFFD; (*aktu&#xFFFD; (*aktu&#xFFFD; (*aktu&#xFFFD; (*aktu&#xFFFD; (*aktu&#xFFFD; (*aktu&#xFFFD; (*aktu&#xFFFD; (*aktu&#xFFFD; (*aktu&#xFFFD; (*aktu&#xFFFD; (*aktu&#xFFFD; (*aktu&#xFFFD; (*aktu&#xFFFD; (*aktu&#xFFFD; (*aktu&#xFFFD; (*aktu&#xFFFD; (*aktu&#xFFFD; (*aktu&#xFFFD; (*aktu&#xFFFD; (*aktu&#xFFFD; (*aktu&#xFFFD; (*aktu&#xFFFD; (*aktu&#xFFFD; (*aktu&#xFFFD; (*aktu&#xFFFD; (*aktu&#xFFFD; (*aktu&#xFFFD; (*aktu&#xFFFD; (*aktu&#xFFFD; (*aktu&#xFFFD; (*aktu&#xFFFD; (*aktu&#xFFFD; (*aktu&#xFFFD; (*aktu&#xFFFD; (*aktu&#xFFFD; (*aktu&#xFFFD; (*aktu&#xFFFD; (*aktu&#xFFFD; (*aktu&#xFFFD; (*aktu&#xFFFD; (*aktu&#xFFFD; (*aktu&#xFFFD; (*aktu&#xFFFD; (*aktu&#xFFFD; (*aktu&#xFFFD; (*aktu&#xFFFD; (*aktu&#xFFFD; (*aktu&#xFFFD; (*aktu&#xFFFD; (*aktu&#xFFFD; (*aktu&#xFFFD; (*aktu&#xFFFD; (*aktu&#xFFFD; (*aktu&#xFFFD; (*aktu&#xFFFD; (*aktu&#xFFFD; (*aktu&#xFFFD; (*aktu&#xFFFD; (*aktu&#xFFFD; (*aktu&#xFFFD; (*aktu&#xFFFD; (*aktu&#xFFFD; (*aktu&#xFFFD; (*aktu&#xFFFD; (*aktu&#xFFFD; (*aktu&#xFFFD; (*aktu&#xFFFD; (*aktu&#xFFFD; (*aktu&#xFFFD; (*aktu&#xFFFD; (*aktu&#xFFFD; (*aktu&#xFFFD; (*aktu&#xFFFD; (*aktu&#xFFFD; (*aktu&#xFFFD; (*aktu&#xFFFD; (*aktu&#xFFFD; (*aktu&#xFFFD; (*aktu&#xFFFD; (*aktu&#xFFFD; (*aktu&#xFFFD; (*aktu&#xFFFD; (*aktu&#xFFFD; (*aktu&#xFFFD; (*aktu&#xFFFD; (*aktu&#xFFFD; (*aktu&#xFFFD; (*aktu&#xFFFD; (*aktu&#xFFFD; (*aktu&#xFFFD; (*aktu&#xFFFD; (*aktu&#xFFFD; (*aktu&#xFFFD; (*aktu&#xFFFD; (*aktu&#xFFFD; (*aktu&#xFFFD; (*aktu&#xFFFD; (*aktu&#xFFFD; (*aktu&#xFFFD; (*aktu&#xFFFD; (*aktu&#xFFFD; (*aktu&#xFFFD; (*aktu&#xFFFD; (*aktu&#xFFFD; (*aktu&#xFFFD; (*aktu&#xFFFD; (*aktu&#xFFFD; (*aktu&#xFFFD; (*aktu&#xFFFD; (*aktu&#xFFFD; (*aktu&#xFFFD; (*aktu&#xFFFD; (*aktu&#xFFFD; (*aktu&#xFFFD; (*aktu&#xFFFD; (*aktu&#xFFFD; (*aktu&#xFFFD; (*aktu&#xFFFD; (*aktu&#xFFFD; (*aktu&#xFFFD; (*aktu&#xFFFD; (*aktu&#xFFFD; (*aktu&#xFFFD; (*aktu&#xFFFD; (*aktu&#xFFFD; (*aktu&#xFFFD; (*aktu&#xFFFD; (*aktu&#xFFFD; (*aktu&#xFFFD; (*aktu&#xFFFD; (*aktu&#xFFFD; (*aktu&#xFFFD; (*aktu&#xFFFD; (*aktu&#xFFFD; (*aktu&#xFFFD; (*aktu&#xFFFD; (*aktu&#xFFFD; (*aktu&#xFFFD; (*aktu&#xFFFD; (*aktu&#xFFFD; (*aktu&#xFFFD; (*aktu&#xFFFD; (*aktu&#xFFFD; (*aktu&#xFFFD; (*aktu&#xFFFD; (*aktu&#xFFFD; (*aktu&#xFFFD; (*aktu&#xFFFD; (*aktu&#xFFFD; (*aktu&#xFFFD; (*aktu&#xFFFD; (*aktu&#xFFFD; (*aktu&#xFFFD; (*aktu&#xFFFD; (*aktu&#xFFFD; (*aktu&#xFFFD; (*aktu&#xFFFD; (*aktu&#xFFFD; (*aktu&#xFFFD; (*aktu&#xFFFD; (*aktu&#xFFFD; (*aktu&#xFFFD; (*aktu&#xFFFD; (*aktu&#xFFFD; (*aktu&#xFFFD; (*aktu&#xFFFD; (*aktu&#xFFFD; (*aktu&#xFFFD; (*aktu&#xFFFD; (*aktu&#xFFFD; (*aktu&#xFFFD; (*aktu&#xFFFD; (*aktu&#xFFFD; (*aktu&#xFFFD; (*aktu&#xFFFD; (*aktu&#xFFFD; (*aktu&#xFFFD; (*aktu&#xFFFD; (*aktu&#xFFFD; (*aktu&#xFFFD; (*aktu&#xFFFD; (*aktu&#xFFFD; (*aktu&#xFFFD; (*aktu&#xFFFD; (*aktu&#xFFFD; (*aktu&#xFFFD; (*aktu&#xFFFD; (*aktu&#xFFFD; (*aktu&#xFFFD; (*aktu&#xFFFD; (*aktu&#xFFFD; (*aktu&#xFFFD; (*aktu&#xFFFD; (*aktu&#xFFFD; (*aktu&#xFFFD; (*aktu&#xFFFD; (*aktu&#xFFFD; (*aktu&#xFFFD; (*aktu&#xFFFD; (*aktu&#xFFFD; (*aktu&#xFFFD; (*aktu&#xFFFD; (*aktu&#xFFFD; (*aktu&#xFFFD; (*aktu&#xFFFD; (*aktu&#xFFFD; (*aktu&#xFFFD; (*aktu&#xFFFD; (*aktu&#xFFFD; (*aktu&#xFFFD; (*aktu&#xFFFD; (*aktu&#xFFFD; (*aktu&#xFFFD; (*aktu&#xFFFD; (*aktu&#xFFFD; (*aktu&#xFFFD; (*aktu&#xFFFD; (*aktu&#xFFFD; (*aktu&#xFFFD; (*aktu&#xFFFD; (*aktu&#xFFFD; (*aktu&#xFFFD; (*aktu&#xFFFD; (*aktu&#xFFFD; (*aktu&#xFFFD; (*aktu&#xFFFD; (*aktu&#xFFFD; (*aktu&#xFFFD; (*aktu&#xFFFD; (*aktu&#xFFFD; (*aktu&#xFFFD; (*aktu&#xFFFD; (*aktu&#xFFFD; (*aktu&#xFFFD; (*aktu&#xFFFD; (*aktu&#xFFFD; (*aktu&#xFFFD; (*aktu&#xFFFD; (*aktu&#xFFFD; (*aktu&#xFFFD; (*aktu&#xFFFD; (*aktu&#xFFFD; (*aktu&#xFFFD; (*aktu&#xFFFD; (*aktu&#xFFFD; (*aktu&#xFFFD; (*aktu&#xFFFD; (*aktu&#xFFFD; (*aktu&#xFFFD; (*aktu&#xFFFD; (*aktu&#xFFFD; (*aktu&#xFFFD; (*aktu&#xFFFD; (*aktu&#xFFFD; (*aktu&#xFFFD; (*aktu&#xFFFD; (*aktu&#xFFFD; (*aktu&#xFFFD; (*aktu&#xFFFD; (*aktu&#xFFFD; (*aktu&#xFFFD; (*aktu&#xFFFD; (*aktu&#xFFFD; (*aktu&#xFFFD; (*aktu&#xFFFD; (*aktu&#xFFFD; (*aktu&#xFFFD; (*aktu&#xFFFD; (*aktu&#xFFFD; (*aktu&#xFFFD; (*aktu&#xFFFD; (*aktu&#xFFFD; (*aktu&#xFFFD; (*aktu&#xFFFD; (*aktu&#xFFFD; (*aktu&#xFFFD; (*aktu&#xFFFD; (*aktu&#xFFFD; (*aktu&#xFFFD; (*aktu&#xFFFD; (*aktu&#xFFFD; (*aktu&#xFFFD; (*aktu&#xFFFD; (*aktu&#xFFFD; (*aktu&#xFFFD; (*aktu&#xFFFD; (*aktu&#xFFFD; (*aktu&#xFFFD; (*aktu&#xFFFD; (*aktu&#xFFFD; (*aktu&#xFFFD; (*aktu&#xFFFD; (*aktu&#xFFFD; (*aktu&#xFFFD; (*aktu&#xFFFD; (*aktu&#xFFFD; (*aktu&#xFFFD; (*aktu&#xFFFD; (*aktu&#xFFFD; (*aktu&#xFFFD; (*aktu&#xFFFD; (*aktu&#xFFFD; (*aktu&#xFFFD; (*aktu&#xFFFD; (*aktu&#xFFFD; (*aktu&#xFFFD; (*aktu&#xFFFD; (*aktu&#xFFFD; (*aktu&#xFFFD; (*aktu&#xFFFD; (*aktu&#xFFFD; (*aktu&#xFFFD; (*aktu&#xFFFD; (*aktu&#xFFFD; (*aktu&#xFFFD; (*aktu&#xFFFD; (*aktu&#xFFFD; (*aktu&#xFFFD; (*aktu&#xFFFD; (*aktu&#xFFFD; (*aktu&#xFFFD; (*aktu&#xFFFD; (*aktu&#xFFFD; (*aktu&#xFFFD; (*aktu&#xFFFD; (*aktu&#xFFFD; (*aktu&#xFFFD; (*aktu&#xFFFD; (*aktu&#xFFFD; (*aktu&#xFFFD; (*aktu&#xFFFD; (*aktu&#xFFFD; (*aktu&#xFFFD; (*aktu&#xFFFD; (*aktu&#xFFFD; (*aktu&#xFFFD; (*aktu&#xFFFD; (*aktu&#xFFFD; (*aktu&#xFFFD; (*aktu&#xFFFD; (*aktu&#xFFFD; (*aktu&#xFFFD; (*aktu&#xFFFD; (*aktu&#xFFFD; (*aktu&#xFFFD; (*aktu&#xFFFD; (*aktu&#xFFFD; (*aktu&#xFFFD; (*aktu&#xFFFD; (*aktu&#xFFFD; (*aktu&#xFFFD; (*aktu&#xFFFD; (*aktu&#xFFFD; (*aktu&#xFFFD; (*aktu&#xFFFD; (*aktu&#xFFFD; (*aktu&#xFFFD; (*aktu&#xFFFD; (*aktu&#xFFFD; (*aktu&#xFFFD; (*aktu&#xFFFD; (*aktu&#xFFFD; (*aktu&#xFFFD; (*aktu&#xFFFD; (*aktu&#xFFFD; (*aktu&#xFFFD; (*aktu&#xFFFD; (*aktu&#xFFFD; (*aktu&#xFFFD; (*aktu&#xFFFD; (*aktu&#xFFFD; (*aktu&#xFFFD; (*aktu&#xFFFD; (*aktu&#xFFFD; (*aktu&#xFFFD; (*aktu&#xFFFD; (*aktu&#xFFFD; (*aktu&#xFFFD; (*aktu&#xFFFD; (*aktu&#xFFFD; (*aktu&#xFFFD; (*aktu&#xFFFD; (*aktu&#xFFFD; (*aktu&#xFFFD; (*aktu&#xFFFD; (*aktu&#xFFFD; (*aktu&#xFFFD; (*aktu&#xFFFD; (*aktu&#xFFFD; (*aktu&#xFFFD; (*aktu&#xFFFD; (*aktu&#xFFFD; (*aktu&#xFFFD; (*aktu&#xFFFD; (*aktu&#xFFFD; (*aktu&#xFFFD; (*aktu&#xFFFD; (*aktu&#xFFFD; (*aktu&#xFFFD; (*aktu&#xFFFD; (*aktu&#xFFFD; (*aktu&#xFFFD; (*aktu&#xFFFD; (*aktu&#xFFFD; (*aktu&#xFFFD; (*aktu&#xFFFD; (*aktu&#xFFFD; (*aktu&#xFFFD; (*aktu&#xFFFD; (*aktu&#xFFFD; (*aktu&#xFFFD; (*aktu&#xFFFD; (*aktu&#xFFFD; (*aktu&#xFFFD; (*aktu&#xFFFD; (*aktu&#xFFFD; (*aktu&#xFFFD; (*aktu&#xFFFD; (*aktu&#xFFFD; (*aktu&#xFFFD; (*aktu&#xFFFD; (*aktu&#xFFFD; (*aktu&#xFFFD; (*aktu&#xFFFD; (*aktu&#xFFFD; (*aktu&#xFFFD; (*aktu&#xFFFD; (*aktu&#xFFFD; (*aktu&#xFFFD; (*aktu&#xFFFD; (*aktu&#xFFFD; (*aktu&#xFFFD; (*aktu&#xFFFD; (*aktu&#xFFFD; (*aktu&#xFFFD; (*aktu&#xFFFD; (*aktu&#xFFFD; (*aktu&#xFFFD; (*aktu&#xFFFD; (*aktu&#xFFFD; (*aktu&#xFFFD; (*aktu&#xFFFD; (*aktu&#xFFFD; (*aktu&#xFFFD; (*aktu&#xFFFD; (*aktu&#xFFFD; (*aktu&#xFFFD; (*aktu&#xFFFD; (*aktu&#xFFFD; (*aktu&#xFFFD; (*aktu&#xFFFD; (*aktu&#xFFFD; (*aktu&#xFFFD; (*aktu&#xFFFD; (*aktu&#xFFFD; (*aktu&#xFFFD; (*aktu&#xFFFD; (*aktu&#xFFFD; (*aktu&#xFFFD; (*aktu&#xFFFD; (*aktu&#xFFFD; (*aktu&#xFFFD; (*aktu&#xFFFD; (*aktu&#xFFFD; (*aktu&#xFFFD; (*aktu&#xFFFD; (*aktu&#xFFFD; (*aktu&#xFFFD; (*aktu&#xFFFD; (*aktu&#xFFFD; (*aktu&#xFFFD; (*aktu&#xFFFD; (*aktu&#xFFFD; (*aktu&#xFFFD; (*aktu&#xFFFD; (*aktu&#xFFFD; (*aktu&#xFFFD; (*aktu&#xFFFD; (*aktu&#xFFFD; (*aktu&#xFFFD; (*aktu&#xFFFD; (*aktu&#xFFFD; (*aktu&#xFFFD; (*aktu&#xFFFD; (*aktu&#xFFFD; (*aktu&#xFFFD; (*aktu&#xFFFD; (*aktu&#xFFFD; (*aktu&#xFFFD; (*aktu&#xFFFD; (*aktu&#xFFFD; (*aktu&#xFFFD; (*aktu&#xFFFD; (*aktu&#xFFFD; (*aktu&#xFFFD; (*aktu&#xFFFD; (*aktu&#xFFFD; (*aktu&#xFFFD; (*aktu&#xFFFD; (*aktu&#xFFFD; (*aktu&#xFFFD; (*aktu&#xFFFD; (*aktu&#xFFFD; (*aktu&#xFFFD; (*aktu&#xFFFD; (*aktu&#xFFFD; (*aktu&#xFFFD; (*aktu&#xFFFD; (*aktu&#xFFFD; (*aktu&#xFFFD; (*aktu&#xFFFD; (*aktu&#xFFFD; (*aktu&#xFFFD; (*aktu&#xFFFD; (*aktu&#xFFFD; (*aktu&#xFFFD; (*aktu&#xFFFD; (*aktu&#xFFFD; (*aktu&#xFFFD; (*aktu&#xFFFD; (*aktu&#xFFFD; (*aktu&#xFFFD; (*aktu&#xFFFD; (*aktu&#xFFFD; (*aktu&#xFFFD; (*aktu&#xFFFD; (*aktu&#xFFFD; (*aktu&#xFFFD; (*aktu&#xFFFD; (*aktu&#xFFFD; (*aktu&#xFFFD; (*aktu&#xFFFD; (*aktu&#xFFFD; (*aktu&#xFFFD; (*aktu&#xFFFD; (*aktu&#xFFFD; (*aktu&#xFFFD; (*aktu&#xFFFD; (*aktu&#xFFFD; (*aktu&#xFFFD; (*aktu&#xFFFD; (*aktu&#xFFFD; (*aktu&#xFFFD; (*aktu&#xFFFD; (*aktu&#xFFFD; (*aktu&#xFFFD; (*aktu&#xFFFD; (*aktu&#xFFFD; (*aktu&#xFFFD; (*aktu&#xFFFD; (*aktu&#xFFFD; (*aktu&#xFFFD; (*aktu&#xFFFD; (*aktu&#xFFFD; (*aktu&#xFFFD; (*aktu&#xFFFD; (*aktu&#xFFFD; (*aktu&#xFFFD; (*aktu&#xFFFD; (*aktu&#xFFFD; (*aktu&#xFFFD; (*aktu&#xFFFD; (*aktu&#xFFFD; (*aktu&#xFFFD; (*aktu&#xFFFD; (*aktu&#xFFFD; (*aktu&#xFFFD; (*aktu&#xFFFD; (*aktu&#xFFFD; (*aktu&#xFFFD; (*aktu&#xFFFD; (*aktu&#xFFFD; (*aktu&#xFFFD; (*aktu&#xFFFD; (*aktu&#xFFFD; (*aktu&#xFFFD; (*aktu&#xFFFD; (*aktu&#xFFFD; (*aktu&#xFFFD; (*aktu&#xFFFD; (*aktu&#xFFFD; (*aktu&#xFFFD; (*aktu&#xFFFD; (*aktu&#xFFFD; (*aktu&#xFFFD; (*aktu&#xFFFD; (*aktu&#xFFFD; (*aktu&#xFFFD; (*aktu&#xFFFD; (*aktu&#xFFFD; (*aktu&#xFFFD; (*aktu&#xFFFD; (*aktu&#xFFFD; (*aktu&#xFFFD; (*aktu&#xFFFD; (*aktu&#xFFFD; (*aktu&#xFFFD; (*aktu&#xFFFD; (*aktu&#xFFFD; (*aktu&#xFFFD; (*aktu&#xFFFD; (*aktu&#xFFFD; (*aktu&#xFFFD; (*aktu&#xFFFD; (*aktu&#xFFFD; (*aktu&#xFFFD; (*aktu&#xFFFD; (*aktu&#xFFFD; (*aktu&#xFFFD; (*aktu&#xFFFD; (*aktu&#xFFFD; (*aktu&#xFFFD; (*aktu&#xFFFD; (*aktu&#xFFFD; (*aktu&#xFFFD; (*aktu&#xFFFD; (*aktu&#xFFFD; (*aktu&#xFFFD; (*aktu&#xFFFD; (*aktu&#xFFFD; (*aktu&#xFFFD; (*aktu&#xFFFD; (*aktu&#xFFFD; (*aktu&#xFFFD; (*aktu&#xFFFD; (*aktu&#xFFFD; (*aktu&#xFFFD; (*aktu&#xFFFD; (*aktu&#xFFFD; (*aktu&#xFFFD; (*aktu&#xFFFD; (*aktu&#xFFFD; (*aktu&#xFFFD; (*aktu&#xFFFD; (*aktu&#xFFFD; (*aktu&#xFFFD; (*aktu&#xFFFD; (*aktu&#xFFFD; (*aktu&#xFFFD; (*aktu&#xFFFD; (*aktu&#xFFFD; (*aktu&#xFFFD; (*aktu&#xFFFD; (*aktu&#xFFFD; (*aktu&#xFFFD; (*aktu&#xFFFD; (*aktu&#xFFFD; (*aktu&#xFFFD; (*aktu&#xFFFD; (*aktu&#xFFFD; (*aktu&#xFFFD; (*aktu&#xFFFD; (*aktu&#xFFFD; (*aktu&#xFFFD; (*aktu&#xFFFD; (*aktu&#xFFFD; (*aktu&#xFFFD; (*aktu&#xFFFD; (*aktu&#xFFFD; (*aktu&#xFFFD; (*aktu&#xFFFD; (*aktu&#xFFFD; (*aktu&#xFFFD; (*aktu&#xFFFD; (*aktu&#xFFFD; (*aktu&#xFFFD; (*aktu&#xFFFD; (*aktu&#xFFFD; (*aktu&#xFFFD; (*aktu&#xFFFD; (*aktu&#xFFFD; (*aktu&#xFFFD; (*aktu&#xFFFD; (*aktu&#xFFFD; (*aktu&#xFFFD; (*aktu&#xFFFD; (*aktu&#xFFFD; (*aktu&#xFFFD; (*aktu&#xFFFD; (*aktu&#xFFFD; (*aktu&#xFFFD; (*aktu&#xFFFD; (*aktu&#xFFFD; (*aktu&#xFFFD; (*aktu&#xFFFD; (*aktu&#xFFFD; (*aktu&#xFFFD; (*aktu&#xFFFD; (*aktu&#xFFFD; (*aktu&#xFFFD; (*aktu&#xFFFD; (*aktu&#xFFFD; (*aktu&#xFFFD; (*aktu&#xFFFD; (*aktu&#xFFFD; (*aktu&#xFFFD; (*aktu&#xFFFD; (*aktu&#xFFFD; (*aktu&#xFFFD; (*aktu&#xFFFD; (*aktu&#xFFFD; (*aktu&#xFFFD; (*aktu&#xFFFD; (*aktu&#xFFFD; (*aktu&#xFFFD; (*aktu&#xFFFD; (*aktu&#xFFFD; (*aktu&#xFFFD; (*aktu&#xFFFD; (*aktu&#xFFFD; (*aktu&#xFFFD; (*aktu&#xFFFD; (*aktu&#xFFFD; (*aktu&#xFFFD; (*aktu&#xFFFD; (*aktu&#xFFFD; (*aktu&#xFFFD; (*aktu&#xFFFD; (*aktu&#xFFFD; (*aktu&#xFFFD; (*aktu&#xFFFD; (*aktu&#xFFFD; (*aktu&#xFFFD; (*aktu&#xFFFD; (*aktu&#xFFFD; (*aktu&#xFFFD; (*aktu&#xFFFD; (*aktu&#xFFFD; (*aktu&#xFFFD; (*aktu&#xFFFD; (*aktu&#xFFFD; (*aktu&#xFFFD; (*aktu&#xFFFD; (*aktu&#xFFFD; (*aktu&#xFFFD; (*aktu&#xFFFD; (*aktu&#xFFFD; (*aktu&#xFFFD; (*aktu&#xFFFD; (*aktu&#xFFFD; (*aktu&#xFFFD; (*aktu&#xFFFD; (*aktu&#xFFFD; (*aktu&#xFFFD; (*aktu&#xFFFD; (*aktu&#xFFFD; (*aktu&#xFFFD; (*aktu&#xFFFD; (*aktu&#xFFFD; (*aktu&#xFFFD; (*aktu&#xFFFD; (*aktu&#xFFFD; (*aktu&#xFFFD; (*aktu&#xFFFD; (*aktu&#xFFFD; (*aktu&#xFFFD; (*aktu&#xFFFD; (*aktu&#xFFFD; (*aktu&#xFFFD; (*aktu&#xFFFD; (*aktu&#xFFFD; (*aktu&#xFFFD; (*aktu&#xFFFD; (*aktu&#xFFFD; (*aktu&#xFFFD; (*aktu&#xFFFD; (*aktu&#xFFFD; (*aktu&#xFFFD; (*aktu&#xFFFD; (*aktu&#xFFFD; (*aktu&#xFFFD; (*aktu&#xFFFD; (*aktu&#xFFFD; (*aktu&#xFFFD; (*aktu&#xFFFD; (*aktu&#xFFFD; (*aktu&#xFFFD; (*aktu&#xFFFD; (*aktu&#xFFFD; (*aktu&#xFFFD; (*aktu&#xFFFD; (*aktu&#xFFFD; (*aktu&#xFFFD; (*aktu&#xFFFD; (*aktu&#xFFFD; (*aktu&#xFFFD; (*aktu&#xFFFD; (*aktu&#xFFFD; (*aktu&#xFFFD; (*aktu&#xFFFD; (*aktu&#xFFFD; (*aktu&#xFFFD; (*aktu&#xFFFD; (*aktu&#xFFFD; (*aktu&#xFFFD; (*aktu&#xFFFD; (*aktu&#xFFFD; (*aktu&#xFFFD; (*aktu&#xFFFD; (*aktu&#xFFFD; (*aktu&#xFFFD; (*aktu&#xFFFD; (*aktu&#xFFFD; (*aktu&#xFFFD; (*aktu&#xFFFD; (*aktu&#xFFFD; (*aktu&#xFFFD; (*aktu&#xFFFD; (*aktu&#xFFFD; (*aktu&#xFFFD; (*aktu&#xFFFD; (*aktu&#xFFFD; (*aktu&#xFFFD; (*aktu&#xFFFD; (*aktu&#xFFFD; (*aktu&#xFFFD; (*aktu&#xFFFD; (*aktu&#xFFFD; (*aktu&#xFFFD; (*aktu&#xFFFD; (*aktu&#xFFFD; (*aktu&#xFFFD; (*aktu&#xFFFD; (*aktu&#xFFFD; (*aktu&#xFFFD; (*aktu&#xFFFD; (*aktu&#xFFFD; (*aktu&#xFFFD; (*aktu&#xFFFD; (*aktu&#xFFFD; (*aktu&#xFFFD; (*aktu&#xFFFD; (*aktu&#xFFFD; (*aktu&#xFFFD; (*aktu&#xFFFD; (*aktu&#xFFFD; (*aktu&#xFFFD; (*aktu&#xFFFD; (*aktu&#xFFFD; (*aktu&#xFFFD; (*aktu&#xFFFD; (*aktu&#xFFFD; (*aktu&#xFFFD; (*aktu&#xFFFD; (*aktu&#xFFFD; (*aktu&#xFFFD; (*aktu&#xFFFD; (*aktu&#xFFFD; (*aktu&#xFFFD; (*aktu&#xFFFD; (*aktu&#xFFFD; (*aktu&#xFFFD; (*aktu&#xFFFD; (*aktu&#xFFFD; (*aktu&#xFFFD; (*aktu&#xFFFD; (*aktu&#xFFFD; (*aktu&#xFFFD; (*aktu&#xFFFD; (*aktu&#xFFFD; (*aktu&#xFFFD; (*aktu&#xFFFD; (*aktu&#xFFFD; (*aktu&#xFFFD; (*aktu&#xFFFD; (*aktu&#xFFFD; (*aktu&#xFFFD; (*aktu&#xFFFD; (*aktu&#xFFFD; (*aktu&#xFFFD; (*aktu&#xFFFD; (*aktu&#xFFFD; (*aktu&#xFFFD; (*aktu&#xFFFD; (*aktu&#xFFFD; (*aktu&#xFFFD; (*aktu&#xFFFD; (*aktu&#xFFFD; (*aktu&#xFFFD; (*aktu&#xFFFD; (*aktu&#xFFFD; (*aktu&#xFFFD; (*aktu&#xFFFD; (*aktu&#xFFFD; (*aktu&#xFFFD; (*aktu&#xFFFD; (*aktu&#xFFFD; (*aktu&#xFFFD; (*aktu&#xFFFD; (*aktu&#xFFFD; (*aktu&#xFFFD; (*aktu&#xFFFD; (*aktu&#xFFFD; (*aktu&#xFFFD; (*aktu&#xFFFD; (*aktu&#xFFFD; (*aktu&#xFFFD; (*aktu&#xFFFD; (*aktu&#xFFFD; (*aktu&#xFFFD; (*aktu&#xFFFD; (*aktu&#xFFFD; (*aktu&#xFFFD; (*aktu&#xFFFD; (*aktu&#xFFFD; (*aktu&#xFFFD; (*aktu&#xFFFD; (*aktu&#xFFFD; (*aktu&#xFFFD; (*aktu&#xFFFD; (*aktu&#xFFFD; (*aktu&#xFFFD; (*aktu&#xFFFD; (*aktu&#xFFFD; (*aktu&#xFFFD; (*aktu&#xFFFD; (*aktu&#xFFFD; (*aktu&#xFFFD; (*aktu&#xFFFD; (*aktu&#xFFFD; (*aktu&#xFFFD; (*aktu&#xFFFD; (*aktu&#xFFFD; (*aktu&#xFFFD; (*aktu&#xFFFD; (*aktu&#xFFFD; (*aktu&#xFFFD; (*aktu&#xFFFD; (*aktu&#xFFFD; (*aktu&#xFFFD; (*aktu&#xFFFD; (*aktu&#xFFFD; (*aktu&#xFFFD; (*aktu&#xFFFD; (*aktu&#xFFFD; (*aktu&#xFFFD; (*aktu&#xFFFD; (*aktu&#xFFFD; (*aktu&#xFFFD; (*aktu&#xFFFD; (*aktu&#xFFFD; (*aktu&#xFFFD; (*aktu&#xFFFD; (*aktu&#xFFFD; (*aktu&#xFFFD; (*aktu&#xFFFD; (*aktu&#xFFFD; (*aktu&#xFFFD; (*aktu&#xFFFD; (*aktu&#xFFFD; (*aktu&#xFFFD; (*aktu&#xFFFD; (*aktu&#xFFFD; (*aktu&#xFFFD; (*aktu&#xFFFD; (*aktu&#xFFFD; (*aktu&#xFFFD; (*aktu&#xFFFD; (*aktu&#xFFFD; (*aktu&#xFFFD; (*aktu&#xFFFD; (*aktu&#xFFFD; (*aktu&#xFFFD; (*aktu&#xFFFD; (*aktu&#xFFFD; (*aktu&#xFFFD; (*aktu&#xFFFD; (*aktu&#xFFFD; (*aktu&#xFFFD; (*aktu&#xFFFD; (*aktu&#xFFFD; (*aktu&#xFFFD; (*aktu&#xFFFD; (*aktu&#xFFFD; (*aktu&#xFFFD; (*aktu&#xFFFD; (*aktu&#xFFFD; (*aktu&#xFFFD; (*aktu&#xFFFD; (*aktu&#xFFFD; (*aktu&#xFFFD; (*aktu&#xFFFD; (*aktu&#xFFFD; (*aktu&#xFFFD; (*aktu&#xFFFD; (*aktu&#xFFFD; (*aktu&#xFFFD; (*aktu&#xFFFD; (*aktu&#xFFFD; (*aktu&#xFFFD; (*aktu&#xFFFD; (*aktu&#xFFFD; (*aktu&#xFFFD; (*aktu&#xFFFD; (*aktu&#xFFFD; (*aktu&#xFFFD; (*aktu&#xFFFD; (*aktu&#xFFFD; (*aktu&#xFFFD; (*aktu&#xFFFD; (*aktu&#xFFFD; (*aktu&#xFFFD; (*aktu&#xFFFD; (*aktu&#xFFFD; (*aktu&#xFFFD; (*aktu&#xFFFD; (*aktu&#xFFFD; (*aktu&#xFFFD; (*aktu&#xFFFD; (*aktu&#xFFFD; (*aktu&#xFFFD; (*aktu&#xFFFD; (*aktu&#xFFFD; (*aktu&#xFFFD; (*aktu&#xFFFD; (*aktu&#xFFFD; (*aktu&#xFFFD; (*aktu&#xFFFD; (*aktu&#xFFFD; (*aktu&#xFFFD; (*aktu&#xFFFD; (*aktu&#xFFFD; (*aktu&#xFFFD; (*aktu&#xFFFD; (*aktu&#xFFFD; (*aktu&#xFFFD; (*aktu&#xFFFD; (*aktu&#xFFFD; (*aktu&#xFFFD; (*aktu&#xFFFD; (*aktu&#xFFFD; (*aktu&#xFFFD; (*aktu&#xFFFD; (*aktu&#xFFFD; (*aktu&#xFFFD; (*aktu&#xFFFD; (*aktu&#xFFFD; (*aktu&#xFFFD; (*aktu&#xFFFD; (*aktu&#xFFFD; (*aktu&#xFFFD; (*aktu&#xFFFD; (*aktu&#xFFFD; (*aktu&#xFFFD; (*aktu&#xFFFD; (*aktu&#xFFFD; (*aktu&#xFFFD; (*aktu&#xFFFD; (*aktu&#xFFFD; (*aktu&#xFFFD; (*aktu&#xFFFD; (*aktu&#xFFFD; (*aktu&#xFFFD; (*aktu&#xFFFD; (*aktu&#xFFFD; (*aktu&#xFFFD; (*aktu&#xFFFD; (*aktu&#xFFFD; (*aktu&#xFFFD; (*aktu&#xFFFD; (*aktu&#xFFFD; (*aktu&#xFFFD; (*aktu&#xFFFD; (*aktu&#xFFFD; (*aktu&#xFFFD; (*aktu&#xFFFD; (*aktu&#xFFFD; (*aktu&#xFFFD; (*aktu&#xFFFD; (*aktu&#xFFFD; (*aktu&#xFFFD; (*aktu&#xFFFD; (*aktu&#xFFFD; (*aktu&#xFFFD; (*aktu&#xFFFD; (*aktu&#xFFFD; (*aktu&#xFFFD; (*aktu&#xFFFD; (*aktu&#xFFFD; (*aktu&#xFFFD; (*aktu&#xFFFD; (*aktu&#xFFFD; (*aktu&#xFFFD; (*aktu&#xFFFD; (*aktu&#xFFFD; (*aktu&#xFFFD; (*aktu&#xFFFD; (*aktu&#xFFFD; (*aktu&#xFFFD; (*aktu&#xFFFD; (*aktu&#xFFFD; (*aktu&#xFFFD; (*aktu&#xFFFD; (*aktu&#xFFFD; (*aktu&#xFFFD; (*aktu&#xFFFD; (*aktu&#xFFFD; (*aktu&#xFFFD; (*aktu&#xFFFD; (*aktu&#xFFFD; (*aktu&#xFFFD; (*aktu&#xFFFD; (*aktu&#xFFFD; (*aktu&#xFFFD; (*aktu&#xFFFD; (*aktu&#xFFFD; (*aktu&#xFFFD; (*aktu&#xFFFD; (*aktu&#xFFFD; (*aktu&#xFFFD; (*aktu&#xFFFD; (*aktu&#xFFFD; (*aktu&#xFFFD; (*aktu&#xFFFD; (*aktu&#xFFFD; (*aktu&#xFFFD; (*aktu&#xFFFD; (*aktu&#xFFFD; (*aktu&#xFFFD; (*aktu&#xFFFD; (*aktu&#xFFFD; (*aktu&#xFFFD; (*aktu&#xFFFD; (*aktu&#xFFFD; (*aktu&#xFFFD; (*aktu&#xFFFD; (*aktu&#xFFFD; (*aktu&#xFFFD; (*aktu&#xFFFD; (*aktu&#xFFFD; (*aktu&#xFFFD; (*aktu&#xFFFD; (*aktu&#xFFFD; (*aktu&#xFFFD; (*aktu&#xFFFD; (*aktu&#xFFFD; (*aktu&#xFFFD; (*aktu&#xFFFD; (*aktu&#xFFFD; (*aktu&#xFFFD; (*aktu&#xFFFD; (*aktu&#xFFFD; (*aktu&#xFFFD; (*aktu&#xFFFD; (*aktu&#xFFFD; (*aktu&#xFFFD; (*aktu&#xFFFD; (*aktu&#xFFFD; (*aktu&#xFFFD; (*aktu&#xFFFD; (*aktu&#xFFFD; (*aktu&#xFFFD; (*aktu&#xFFFD; (*aktu&#xFFFD; (*aktu&#xFFFD; (*aktu&#xFFFD; (*aktu&#xFFFD; (*aktu&#xFFFD; (*aktu&#xFFFD; (*aktu&#xFFFD; (*aktu&#xFFFD; (*aktu&#xFFFD; (*aktu&#xFFFD; (*aktu&#xFFFD; (*aktu&#xFFFD; (*aktu&#xFFFD; (*aktu&#xFFFD; (*aktu&#xFFFD; (*aktu&#xFFFD; (*aktu&#xFFFD; (*aktu&#xFFFD; (*aktu&#xFFFD; (*aktu&#xFFFD; (*aktu&#xFFFD; (*aktu&#xFFFD; (*aktu&#xFFFD; (*aktu&#xFFFD; (*aktu&#xFFFD; (*aktu&#xFFFD; (*aktu&#xFFFD; (*aktu&#xFFFD; (*aktu&#xFFFD; (*aktu&#xFFFD; (*aktu&#xFFFD; (*aktu&#xFFFD; (*aktu&#xFFFD; (*aktu&#xFFFD; (*aktu&#xFFFD; (*aktu&#xFFFD; (*aktu&#xFFFD; (*aktu&#xFFFD; (*aktu&#xFFFD; (*aktu&#xFFFD; (*aktu&#xFFFD; (*aktu&#xFFFD; (*aktu&#xFFFD; (*aktu&#xFFFD; (*aktu&#xFFFD; (*aktu&#xFFFD; (*aktu&#xFFFD; (*aktu&#xFFFD; (*aktu&#xFFFD; (*aktu&#xFFFD; (*aktu&#xFFFD; (*aktu&#xFFFD; (*aktu&#xFFFD; (*aktu&#xFFFD; (*aktu&#xFFFD; (*aktu&#xFFFD; (*aktu&#xFFFD; (*aktu&#xFFFD; (*aktu&#xFFFD; (*aktu&#xFFFD; (*aktu&#xFFFD; (*aktu&#xFFFD; (*aktu&#xFFFD; (*aktu&#xFFFD; (*aktu&#xFFFD; (*aktu&#xFFFD; (*aktu&#xFFFD; (*aktu&#xFFFD; (*aktu&#xFFFD; (*aktu&#xFFFD; (*aktu&#xFFFD; (*aktu&#xFFFD; (*aktu&#xFFFD; (*aktu&#xFFFD; (*aktu&#xFFFD; (*aktu&#xFFFD; (*aktu&#xFFFD; (*aktu&#xFFFD; (*aktu&#xFFFD; (*aktu&#xFFFD; (*aktu&#xFFFD; (*aktu&#xFFFD; (*aktu&#xFFFD; (*aktu&#xFFFD; (*aktu&#xFFFD; (*aktu&#xFFFD; (*aktu&#xFFFD; (*aktu&#xFFFD; (*aktu&#xFFFD; (*aktu&#xFFFD; (*aktu&#xFFFD; (*aktu&#xFFFD; (*aktu&#xFFFD; (*aktu&#xFFFD; (*aktu&#xFFFD; (*aktu&#xFFFD; (*aktu&#xFFFD; (*aktu&#xFFFD; (*aktu&#xFFFD; (*aktu&#xFFFD; (*aktu&#xFFFD; (*aktu&#xFFFD; (*aktu&#xFFFD; (*aktu&#xFFFD; (*aktu&#xFFFD; (*aktu&#xFFFD; (*aktu&#xFFFD; (*aktu&#xFFFD; (*aktu&#xFFFD; (*aktu&#xFFFD; (*aktu&#xFFFD; (*aktu&#xFFFD; (*aktu&#xFFFD; (*aktu&#xFFFD; (*aktu&#xFFFD; (*aktu&#xFFFD; (*aktu&#xFFFD; (*aktu&#xFFFD; (*aktu&#xFFFD; (*aktu&#xFFFD; (*aktu&#xFFFD; (*aktu&#xFFFD; (*aktu&#xFFFD; (*aktu&#xFFFD; (*aktu&#xFFFD; (*aktu&#xFFFD; (*aktu&#xFFFD; (*aktu&#xFFFD; (*aktu&#xFFFD; (*aktu&#xFFFD; (*aktu&#xFFFD; (*aktu&#xFFFD; (*aktu&#xFFFD; (*aktu&#xFFFD; (*aktu&#xFFFD; (*aktu&#xFFFD; (*aktu&#xFFFD; (*aktu&#xFFFD; (*aktu&#xFFFD; (*aktu&#xFFFD; (*aktu&#xFFFD; (*aktu&#xFFFD; (*aktu&#xFFFD; (*aktu&#xFFFD; (*aktu&#xFFFD; (*aktu&#xFFFD; (*aktu&#xFFFD; (*aktu&#xFFFD; (*aktu&#xFFFD; (*aktu&#xFFFD; (*aktu&#xFFFD; (*aktu&#xFFFD; (*aktu&#xFFFD; (*aktu&#xFFFD; (*aktu&#xFFFD; (*aktu&#xFFFD; (*aktu&#xFFFD; (*aktu&#xFFFD; (*aktu&#xFFFD; (*aktu&#xFFFD; (*aktu&#xFFFD; (*aktu&#xFFFD; (*aktu&#xFFFD; (*aktu&#xFFFD; (*aktu&#xFFFD; (*aktu&#xFFFD; (*aktu&#xFFFD; (*aktu&#xFFFD; (*aktu&#xFFFD; (*aktu&#xFFFD; (*aktu&#xFFFD; (*aktu&#xFFFD; (*aktu&#xFFFD; (*aktu&#xFFFD; (*aktu&#xFFFD; (*aktu&#xFFFD; (*aktu&#xFFFD; (*aktu&#xFFFD; (*aktu&#xFFFD; (*aktu&#xFFFD; (*aktu&#xFFFD; (*aktu&#xFFFD; (*aktu&#xFFFD; (*aktu&#xFFFD; (*aktu&#xFFFD; (*aktu&#xFFFD; (*aktu&#xFFFD; (*aktu&#xFFFD; (*aktu&#xFFFD; (*aktu&#xFFFD; (*aktu&#xFFFD; (*aktu&#xFFFD; (*aktu&#xFFFD; (*aktu&#xFFFD; (*aktu&#xFFFD; (*aktu&#xFFFD; (*aktu&#xFFFD; (*aktu&#xFFFD; (*aktu&#xFFFD; (*aktu&#xFFFD; (*aktu&#xFFFD; (*aktu&#xFFFD; (*aktu&#xFFFD; (*aktu&#xFFFD; (*aktu&#xFFFD; (*aktu&#xFFFD; (*aktu&#xFFFD; (*aktu&#xFFFD; (*aktu&#xFFFD; (*aktu&#xFFFD; (*aktu&#xFFFD; (*aktu&#xFFFD; (*aktu&#xFFFD; (*aktu&#xFFFD; (*aktu&#xFFFD; (*aktu&#xFFFD; (*aktu&#xFFFD; (*aktu&#xFFFD; (*aktu&#xFFFD; (*aktu&#xFFFD; (*aktu&#xFFFD; (*aktu&#xFFFD; (*aktu&#xFFFD; (*aktu&#xFFFD; (*aktu&#xFFFD; (*aktu&#xFFFD; (*aktu&#xFFFD; (*aktu&#xFFFD; (*aktu&#xFFFD; (*aktu&#xFFFD; (*aktu&#xFFFD; (*aktu&#xFFFD; (*aktu&#xFFFD; (*aktu&#xFFFD; (*aktu&#xFFFD; (*aktu&#xFFFD; (*aktu&#xFFFD; (*aktu&#xFFFD; (*aktu&#xFFFD; (*aktu&#xFFFD; (*aktu&#xFFFD; (*aktu&#xFFFD; (*aktu&#xFFFD; (*aktu&#xFFFD; (*aktu&#xFFFD; (*aktu&#xFFFD; (*aktu&#xFFFD; (*aktu&#xFFFD; (*aktu&#xFFFD; (*aktu&#xFFFD; (*aktu&#xFFFD; (*aktu&#xFFFD; (*aktu&#xFFFD; (*aktu&#xFFFD; (*aktu&#xFFFD; (*aktu&#xFFFD; (*aktu&#xFFFD; (*aktu&#xFFFD; (*aktu&#xFFFD; (*aktu&#xFFFD; (*aktu&#xFFFD; (*aktu&#xFFFD; (*aktu&#xFFFD; (*aktu&#xFFFD; (*aktu&#xFFFD; (*aktu&#xFFFD; (*aktu&#xFFFD; (*aktu&#xFFFD; (*aktu&#xFFFD; (*aktu&#xFFFD; (*aktu&#xFFFD; (*aktu&#xFFFD; (*aktu&#xFFFD; (*aktu&#xFFFD; (*aktu&#xFFFD; (*aktu&#xFFFD; (*aktu&#xFFFD; (*aktu&#xFFFD; (*aktu&#xFFFD; (*aktu&#xFFFD; (*aktu&#xFFFD; (*aktu&#xFFFD; (*aktu&#xFFFD; (*aktu&#xFFFD; (*aktu&#xFFFD; (*aktu&#xFFFD; (*aktu&#xFFFD; (*aktu&#xFFFD; (*aktu&#xFFFD; (*aktu&#xFFFD; (*aktu&#xFFFD; (*aktu&#xFFFD; (*aktu&#xFFFD; (*aktu&#xFFFD; (*aktu&#xFFFD; (*aktu&#xFFFD; (*aktu&#xFFFD; (*aktu&#xFFFD; (*aktu&#xFFFD; (*aktu&#xFFFD; (*aktu&#xFFFD; (*aktu&#xFFFD; (*aktu&#xFFFD; (*aktu&#xFFFD; (*aktu&#xFFFD; (*aktu&#xFFFD; (*aktu&#xFFFD; (*aktu&#xFFFD; (*aktu&#xFFFD; (*aktu&#xFFFD; (*aktu&#xFFFD; (*aktu&#xFFFD; (*aktu&#xFFFD; (*aktu&#xFFFD; (*aktu&#xFFFD; (*aktu&#xFFFD; (*aktu&#xFFFD; (*aktu&#xFFFD; (*aktu&#xFFFD; (*aktu&#xFFFD; (*aktu&#xFFFD; (*aktu&#xFFFD; (*aktu&#xFFFD; (*aktu&#xFFFD; (*aktu&#xFFFD; (*aktu&#xFFFD; (*aktu&#xFFFD; (*aktu&#xFFFD; (*aktu&#xFFFD; (*aktu&#xFFFD; (*aktu&#xFFFD; (*aktu&#xFFFD; (*aktu&#xFFFD; (*aktu&#xFFFD; (*aktu&#xFFFD; (*aktu&#xFFFD; (*aktu&#xFFFD; (*aktu&#xFFFD; (*aktu&#xFFFD; (*aktu&#xFFFD; (*aktu&#xFFFD; (*aktu&#xFFFD; (*aktu&#xFFFD; (*aktu&#xFFFD; (*aktu&#xFFFD; (*aktu&#xFFFD; (*aktu&#xFFFD; (*aktu&#xFFFD; (*aktu&#xFFFD; (*aktu&#xFFFD; (*aktu&#xFFFD; (*aktu&#xFFFD; (*aktu&#xFFFD; (*aktu&#xFFFD; (*aktu&#xFFFD; (*aktu&#xFFFD; (*aktu&#xFFFD; (*aktu&#xFFFD; (*aktu&#xFFFD; (*aktu&#xFFFD; (*aktu&#xFFFD; (*aktu&#xFFFD; (*aktu&#xFFFD; (*aktu&#xFFFD; (*aktu&#xFFFD; (*aktu&#xFFFD; (*aktu&#xFFFD; (*aktu&#xFFFD; (*aktu&#xFFFD; (*aktu&#xFFFD; (*aktu&#xFFFD; (*aktu&#xFFFD; (*aktu&#xFFFD; (*aktu&#xFFFD; (*aktu&#xFFFD; (*aktu&#xFFFD; (*aktu&#xFFFD; (*aktu&#xFFFD; (*aktu&#xFFFD; (*aktu&#xFFFD; (*aktu&#xFFFD; (*aktu&#xFFFD; (*aktu&#xFFFD; (*aktu&#xFFFD; (*aktu&#xFFFD; (*aktu&#xFFFD; (*aktu&#xFFFD; (*aktu&#xFFFD; (*aktu&#xFFFD; (*aktu&#xFFFD; (*aktu&#xFFFD; (*aktu&#xFFFD; (*aktu&#xFFFD; (*aktu&#xFFFD; (*aktu&#xFFFD; (*aktu&#xFFFD; (*aktu&#xFFFD; (*aktu&#xFFFD; (*aktu&#xFFFD; (*aktu&#xFFFD; (*aktu&#xFFFD; (*aktu&#xFFFD; (*aktu&#xFFFD; (*aktu&#xFFFD; (*aktu&#xFFFD; (*aktu&#xFFFD; (*aktu&#xFFFD; (*aktu&#xFFFD; (*aktu&#xFFFD; (*aktu&#xFFFD; (*aktu&#xFFFD; (*aktu&#xFFFD; (*aktu&#xFFFD; (*aktu&#xFFFD; (*aktu&#xFFFD; (*aktu&#xFFFD; (*aktu&#xFFFD; (*aktu&#xFFFD; (*aktu&#xFFFD; (*aktu&#xFFFD; (*aktu&#xFFFD; (*aktu&#xFFFD; (*aktu&#xFFFD; (*aktu&#xFFFD; (*aktu&#xFFFD; (*aktu&#xFFFD; (*aktu&#xFFFD; (*aktu&#xFFFD; (*aktu&#xFFFD; (*aktu&#xFFFD; (*aktu&#xFFFD; (*aktu&#xFFFD; (*aktu&#xFFFD; (*aktu&#xFFFD; (*aktu&#xFFFD; (*aktu&#xFFFD; (*aktu&#xFFFD; (*aktu&#xFFFD; (*aktu&#xFFFD; (*aktu&#xFFFD; (*aktu&#xFFFD; (*aktu&#xFFFD; (*aktu&#xFFFD; (*aktu&#xFFFD; (*aktu&#xFFFD; (*aktu&#xFFFD; (*aktu&#xFFFD; (*aktu&#xFFFD; (*aktu&#xFFFD; (*aktu&#xFFFD; (*aktu&#xFFFD; (*aktu&#xFFFD; (*aktu&#xFFFD; (*aktu&#xFFFD; (*aktu&#xFFFD; (*aktu&#xFFFD; (*aktu&#xFFFD; (*aktu&#xFFFD; (*aktu&#xFFFD; (*aktu&#xFFFD; (*aktu&#xFFFD; (*aktu&#xFFFD; (*aktu&#xFFFD; (*aktu&#xFFFD; (*aktu&#xFFFD; (*aktu&#xFFFD; (*aktu&#xFFFD; (*aktu&#xFFFD; (*aktu&#xFFFD; (*aktu&#xFFFD; (*aktu&#xFFFD; (*aktu&#xFFFD; (*aktu&#xFFFD; (*aktu&#xFFFD; (*aktu&#xFFFD; (*aktu&#xFFFD; (*aktu&#xFFFD; (*aktu&#xFFFD; (*aktu&#xFFFD; (*aktu&#xFFFD; (*aktu&#xFFFD; (*aktu&#xFFFD; (*aktu&#xFFFD; (*aktu&#xFFFD; (*aktu&#xFFFD; (*aktu&#xFFFD; (*aktu&#xFFFD; (*aktu&#xFFFD; (*aktu&#xFFFD; (*aktu&#xFFFD; (*aktu&#xFFFD; (*aktu&#xFFFD; (*aktu&#xFFFD; (*aktu&#xFFFD; (*aktu&#xFFFD; (*aktu&#xFFFD; (*aktu&#xFFFD; (*aktu&#xFFFD; (*aktu&#xFFFD; (*aktu&#xFFFD; (*aktu&#xFFFD; (*aktu&#xFFFD; (*aktu&#xFFFD; (*aktu&#xFFFD; (*aktu&#xFFFD; (*aktu&#xFFFD; (*aktu&#xFFFD; (*aktu&#xFFFD; (*aktu&#xFFFD; (*aktu&#xFFFD; (*aktu&#xFFFD; (*aktu&#xFFFD; (*aktu&#xFFFD; (*aktu&#xFFFD; (*aktu&#xFFFD; (*aktu&#xFFFD; (*aktu&#xFFFD; (*aktu&#xFFFD; (*aktu&#xFFFD; (*aktu&#xFFFD; (*aktu&#xFFFD; (*aktu&#xFFFD; (*aktu&#xFFFD; (*aktu&#xFFFD; (*aktu&#xFFFD; (*aktu&#xFFFD; (*aktu&#xFFFD; (*aktu&#xFFFD; (*aktu&#xFFFD; (*aktu&#xFFFD; (*aktu&#xFFFD; (*aktu&#xFFFD; (*aktu&#xFFFD; (*aktu&#xFFFD; (*aktu&#xFFFD; (*aktu&#xFFFD; (*aktu&#xFFFD; (*aktu&#xFFFD; (*aktu&#xFFFD; (*aktu&#xFFFD; (*aktu&#xFFFD; (*aktu&#xFFFD; (*aktu&#xFFFD; (*aktu&#xFFFD; (*aktu&#xFFFD; (*aktu&#xFFFD; (*aktu&#xFFFD; (*aktu&#xFFFD; (*aktu&#xFFFD; (*aktu&#xFFFD; (*aktu&#xFFFD; (*aktu&#xFFFD; (*aktu&#xFFFD; (*aktu&#xFFFD; (*aktu&#xFFFD; (*aktu&#xFFFD; (*aktu&#xFFFD; (*aktu&#xFFFD; (*aktu&#xFFFD; (*aktu&#xFFFD; (*aktu&#xFFFD; (*aktu&#xFFFD; (*aktu&#xFFFD; (*aktu&#xFFFD; (*aktu&#xFFFD; (*aktu&#xFFFD; (*aktu&#xFFFD; (*aktu&#xFFFD; (*aktu&#xFFFD; (*aktu&#xFFFD; (*aktu&#xFFFD; (*aktu&#xFFFD; (*aktu&#xFFFD; (*aktu&#xFFFD; (*aktu&#xFFFD; (*aktu&#xFFFD; (*aktu&#xFFFD; (*aktu&#xFFFD; (*aktu&#xFFFD; (*aktu&#xFFFD; (*aktu&#xFFFD; (*aktu&#xFFFD; (*aktu&#xFFFD; (*aktu&#xFFFD; (*aktu&#xFFFD; (*aktu&#xFFFD; (*aktu&#xFFFD; (*aktu&#xFFFD; (*aktu&#xFFFD; (*aktu&#xFFFD; (*aktu&#xFFFD; (*aktu&#xFFFD; (*aktu&#xFFFD; (*aktu&#xFFFD; (*aktu&#xFFFD; (*aktu&#xFFFD; (*aktu&#xFFFD; (*aktu&#xFFFD; (*aktu&#xFFFD; (*aktu&#xFFFD; (*aktu&#xFFFD; (*aktu&#xFFFD; (*aktu&#xFFFD; (*aktu&#xFFFD; (*aktu&#xFFFD; (*aktu&#xFFFD; (*aktu&#xFFFD; (*aktu&#xFFFD; (*aktu&#xFFFD; (*aktu&#xFFFD; (*aktu&#xFFFD; (*aktu&#xFFFD; (*aktu&#xFFFD; (*aktu&#xFFFD; (*aktu&#xFFFD; (*aktu&#xFFFD; (*aktu&#xFFFD; (*aktu&#xFFFD; (*aktu&#xFFFD; (*aktu&#xFFFD; (*aktu&#xFFFD; (*aktu&#xFFFD; (*aktu&#xFFFD; (*aktu&#xFFFD; (*aktu&#xFFFD; (*aktu&#xFFFD; (*aktu&#xFFFD; (*aktu&#xFFFD; (*aktu&#xFFFD; (*aktu&#xFFFD; (*aktu&#xFFFD; (*aktu&#xFFFD; (*aktu&#xFFFD; (*aktu&#xFFFD; (*aktu&#xFFFD; (*aktu&#xFFFD; (*aktu&#xFFFD; (*aktu&#xFFFD; (*aktu&#xFFFD; (*aktu&#xFFFD; (*aktu&#xFFFD; (*aktu&#xFFFD; (*aktu&#xFFFD; (*aktu&#xFFFD; (*aktu&#xFFFD; (*aktu&#xFFFD; (*aktu&#xFFFD; (*aktu&#xFFFD; (*aktu&#xFFFD; (*aktu&#xFFFD; (*aktu&#xFFFD; (*aktu&#xFFFD; (*aktu&#xFFFD; (*aktu&#xFFFD; (*aktu&#xFFFD; (*aktu&#xFFFD; (*aktu&#xFFFD; (*aktu&#xFFFD; (*aktu&#xFFFD; (*aktu&#xFFFD; (*aktu&#xFFFD; (*aktu&#xFFFD; (*aktu&#xFFFD; (*aktu&#xFFFD; (*aktu&#xFFFD; (*aktu&#xFFFD; (*aktu&#xFFFD; (*aktu&#xFFFD; (*aktu&#xFFFD; (*aktu&#xFFFD; (*aktu&#xFFFD; (*aktu&#xFFFD; (*aktu&#xFFFD; (*aktu&#xFFFD; (*aktu&#xFFFD; (*aktu&#xFFFD; (*aktu&#xFFFD; (*aktu&#xFFFD; (*aktu&#xFFFD; (*aktu&#xFFFD; (*aktu&#xFFFD; (*aktu&#xFFFD; (*aktu&#xFFFD; (*aktu&#xFFFD; (*aktu&#xFFFD; (*aktu&#xFFFD; (*aktu&#xFFFD; (*aktu&#xFFFD; (*aktu&#xFFFD; (*aktu&#xFFFD; (*aktu&#xFFFD; (*aktu&#xFFFD; (*aktu&#xFFFD; (*aktu&#xFFFD; (*aktu&#xFFFD; (*aktu&#xFFFD; (*aktu&#xFFFD; (*aktu&#xFFFD; (*aktu&#xFFFD; (*aktu&#xFFFD; (*aktu&#xFFFD; (*aktu&#xFFFD; (*aktu&#xFFFD; (*aktu&#xFFFD; (*aktu&#xFFFD; (*aktu&#xFFFD; (*aktu&#xFFFD; (*aktu&#xFFFD; (*aktu&#xFFFD; (*aktu&#xFFFD; (*aktu&#xFFFD; (*aktu&#xFFFD; (*aktu&#xFFFD; (*aktu&#xFFFD; (*aktu&#xFFFD; (*aktu&#xFFFD; (*aktu&#xFFFD; (*aktu&#xFFFD; (*aktu&#xFFFD; (*aktu&#xFFFD; (*aktu&#xFFFD; (*aktu&#xFFFD; (*aktu&#xFFFD; (*aktu&#xFFFD; (*aktu&#xFFFD; (*aktu&#xFFFD; (*aktu&#xFFFD; (*aktu&#xFFFD; (*aktu&#xFFFD; (*aktu&#xFFFD; (*aktu&#xFFFD; (*aktu&#xFFFD; (*aktu&#xFFFD; (*aktu&#xFFFD; (*aktu&#xFFFD; (*aktu&#xFFFD; (*aktu&#xFFFD; (*aktu&#xFFFD; (*aktu&#xFFFD; (*aktu&#xFFFD; (*aktu&#xFFFD; (*aktu&#xFFFD; (*aktu&#xFFFD; (*aktu&#xFFFD; (*aktu&#xFFFD; (*aktu&#xFFFD; (*aktu&#xFFFD; (*aktu&#xFFFD; (*aktu&#xFFFD; (*aktu&#xFFFD; (*aktu&#xFFFD; (*aktu&#xFFFD; (*aktu&#xFFFD; (*aktu&#xFFFD; (*aktu&#xFFFD; (*aktu&#xFFFD; (*aktu&#xFFFD; (*aktu&#xFFFD; (*aktu&#xFFFD; (*aktu&#xFFFD; (*aktu&#xFFFD; (*aktu&#xFFFD; (*aktu&#xFFFD; (*aktu&#xFFFD; (*aktu&#xFFFD; (*aktu&#xFFFD; (*aktu&#xFFFD; (*aktu&#xFFFD; (*aktu&#xFFFD; (*aktu&#xFFFD; (*aktu&#xFFFD; (*aktu&#xFFFD; (*aktu&#xFFFD; (*aktu&#xFFFD; (*aktu&#xFFFD; (*aktu&#xFFFD; (*aktu&#xFFFD; (*aktu&#xFFFD; (*aktu&#xFFFD; (*aktu&#xFFFD; (*aktu&#xFFFD; (*aktu&#xFFFD; (*aktu&#xFFFD; (*aktu&#xFFFD; (*aktu&#xFFFD; (*aktu&#xFFFD; (*aktu&#xFFFD; (*aktu&#xFFFD; (*aktu&#xFFFD; (*aktu&#xFFFD; (*aktu&#xFFFD; (*aktu&#xFFFD; (*aktu&#xFFFD; (*aktu&#xFFFD; (*aktu&#xFFFD; (*aktu&#xFFFD; (*aktu&#xFFFD; (*aktu&#xFFFD; (*aktu&#xFFFD; (*aktu&#xFFFD; (*aktu&#xFFFD; (*aktu&#xFFFD; (*aktu&#xFFFD; (*aktu&#xFFFD; (*aktu&#xFFFD; (*aktu&#xFFFD; (*aktu&#xFFFD; (*aktu&#xFFFD; (*aktu&#xFFFD; (*aktu&#xFFFD; (*aktu&#xFFFD; (*aktu&#xFFFD; (*aktu&#xFFFD; (*aktu&#xFFFD; (*aktu&#xFFFD; (*aktu&#xFFFD; (*aktu&#xFFFD; (*aktu&#xFFFD; (*aktu&#xFFFD; (*aktu&#xFFFD; (*aktu&#xFFFD; (*aktu&#xFFFD; (*aktu&#xFFFD; (*aktu&#xFFFD; (*aktu&#xFFFD; (*aktu&#xFFFD; (*aktu&#xFFFD; (*aktu&#xFFFD; (*aktu&#xFFFD; (*aktu&#xFFFD; (*aktu&#xFFFD; (*aktu&#xFFFD; (*aktu&#xFFFD; (*aktu&#xFFFD; (*aktu&#xFFFD; (*aktu&#xFFFD; (*aktu&#xFFFD; (*aktu&#xFFFD; (*aktu&#xFFFD; (*aktu&#xFFFD; (*aktu&#xFFFD; (*aktu&#xFFFD; (*aktu&#xFFFD; (*aktu&#xFFFD; (*aktu&#xFFFD; (*aktu&#xFFFD; (*aktu&#xFFFD; (*aktu&#xFFFD; (*aktu&#xFFFD; (*aktu&#xFFFD; (*aktu&#xFFFD; (*aktu&#xFFFD; (*aktu&#xFFFD; (*aktu&#xFFFD; (*aktu&#xFFFD; (*aktu&#xFFFD; (*aktu&#xFFFD; (*aktu&#xFFFD; (*aktu&#xFFFD; (*aktu&#xFFFD; (*aktu&#xFFFD; (*aktu&#xFFFD; (*aktu&#xFFFD; (*aktu&#xFFFD; (*aktu&#xFFFD; (*aktu&#xFFFD; (*aktu&#xFFFD; (*aktu&#xFFFD; (*aktu&#xFFFD; (*aktu&#xFFFD; (*aktu&#xFFFD; (*aktu&#xFFFD; (*aktu&#xFFFD; (*aktu&#xFFFD; (*aktu&#xFFFD; (*aktu&#xFFFD; (*aktu&#xFFFD; (*aktu&#xFFFD; (*aktu&#xFFFD; (*aktu&#xFFFD; (*aktu&#xFFFD; (*aktu&#xFFFD; (*aktu&#xFFFD; (*aktu&#xFFFD; (*aktu&#xFFFD; (*aktu&#xFFFD; (*aktu&#xFFFD; (*aktu&#xFFFD; (*aktu&#xFFFD; (*aktu&#xFFFD; (*aktu&#xFFFD; (*aktu&#xFFFD; (*aktu&#xFFFD; (*aktu&#xFFFD; (*aktu&#xFFFD; (*aktu&#xFFFD; (*aktu&#xFFFD; (*aktu&#xFFFD; (*aktu&#xFFFD; (*aktu&#xFFFD; (*aktu&#xFFFD; (*aktu&#xFFFD; (*aktu&#xFFFD; (*aktu&#xFFFD; (*aktu&#xFFFD; (*aktu&#xFFFD; (*aktu&#xFFFD; (*aktu&#xFFFD; (*aktu&#xFFFD; (*aktu&#xFFFD; (*aktu&#xFFFD; (*aktu&#xFFFD; (*aktu&#xFFFD; (*aktu&#xFFFD; (*aktu&#xFFFD; (*aktu&#xFFFD; (*aktu&#xFFFD; (*aktu&#xFFFD; (*aktu&#xFFFD; (*aktu&#xFFFD; (*aktu&#xFFFD; (*aktu&#xFFFD; (*aktu&#xFFFD; (*aktu&#xFFFD; (*aktu&#xFFFD; (*aktu&#xFFFD; (*aktu&#xFFFD; (*aktu&#xFFFD; (*aktu&#xFFFD; (*aktu&#xFFFD; (*aktu&#xFFFD; (*aktu&#xFFFD; (*aktu&#xFFFD; (*aktu&#xFFFD; (*aktu&#xFFFD; (*aktu&#xFFFD; (*aktu&#xFFFD; (*aktu&#xFFFD; (*aktu&#xFFFD; (*aktu&#xFFFD; (*aktu&#xFFFD; (*aktu&#xFFFD; (*aktu&#xFFFD; (*aktu&#xFFFD; (*aktu&#xFFFD; (*aktu&#xFFFD; (*aktu&#xFFFD; (*aktu&#xFFFD; (*aktu&#xFFFD; (*aktu&#xFFFD; (*aktu&#xFFFD; (*aktu&#xFFFD; (*aktu&#xFFFD; (*aktu&#xFFFD; (*aktu&#xFFFD; (*aktu&#xFFFD; (*aktu&#xFFFD; (*aktu&#xFFFD; (*aktu&#xFFFD; (*aktu&#xFFFD; (*aktu&#xFFFD; (*aktu&#xFFFD; (*aktu&#xFFFD; (*aktu&#xFFFD; (*aktu&#xFFFD; (*aktu&#xFFFD; (*aktu&#xFFFD; (*aktu&#xFFFD; (*aktu&#xFFFD; (*aktu&#xFFFD; (*aktu&#xFFFD; (*aktu&#xFFFD; (*aktu&#xFFFD; (*aktu&#xFFFD; (*aktu&#xFFFD; (*aktu&#xFFFD; (*aktu&#xFFFD; (*aktu&#xFFFD; (*aktu&#xFFFD; (*aktu&#xFFFD; (*aktu&#xFFFD; (*aktu&#xFFFD; (*aktu&#xFFFD; (*aktu&#xFFFD; (*aktu&#xFFFD; (*aktu&#xFFFD; (*aktu&#xFFFD; (*aktu&#xFFFD; (*aktu&#xFFFD; (*aktu&#xFFFD; (*aktu&#xFFFD; (*aktu&#xFFFD; (*aktu&#xFFFD; (*aktu&#xFFFD; (*aktu&#xFFFD; (*aktu&#xFFFD; (*aktu&#xFFFD; (*aktu&#xFFFD; (*aktu&#xFFFD; (*aktu&#xFFFD; (*aktu&#xFFFD; (*aktu&#xFFFD; (*aktu&#xFFFD; (*aktu&#xFFFD; (*aktu&#xFFFD; (*aktu&#xFFFD; (*aktu&#xFFFD; (*aktu&#xFFFD; (*aktu&#xFFFD; (*aktu&#xFFFD; (*aktu&#xFFFD; (*aktu&#xFFFD; (*aktu&#xFFFD; (*aktu&#xFFFD; (*aktu&#xFFFD; (*aktu&#xFFFD; (*aktu&#xFFFD; (*aktu&#xFFFD; (*aktu&#xFFFD; (*aktu&#xFFFD; (*aktu&#xFFFD; (*aktu&#xFFFD; (*aktu&#xFFFD; (*aktu&#xFFFD; (*aktu&#xFFFD; (*aktu&#xFFFD; (*aktu&#xFFFD; (*aktu&#xFFFD; (*aktu&#xFFFD; (*aktu&#xFFFD; (*aktu&#xFFFD; (*aktu&#xFFFD; (*aktu&#xFFFD; (*aktu&#xFFFD; (*aktu&#xFFFD; (*aktu&#xFFFD; (*aktu&#xFFFD; (*aktu&#xFFFD; (*aktu&#xFFFD; (*aktu&#xFFFD; (*aktu&#xFFFD; (*aktu&#xFFFD; (*aktu&#xFFFD; (*aktu&#xFFFD; (*aktu&#xFFFD; (*aktu&#xFFFD; (*aktu&#xFFFD; (*aktu&#xFFFD; (*aktu&#xFFFD; (*aktu&#xFFFD; (*aktu&#xFFFD; (*aktu&#xFFFD; (*aktu&#xFFFD; (*aktu&#xFFFD; (*aktu&#xFFFD; (*aktu&#xFFFD; (*aktu&#xFFFD; (*aktu&#xFFFD; (*aktu&#xFFFD; (*aktu&#xFFFD; (*aktu&#xFFFD; (*aktu&#xFFFD; (*aktu&#xFFFD; (*aktu&#xFFFD; (*aktu&#xFFFD; (*aktu&#xFFFD; (*aktu&#xFFFD; (*aktu&#xFFFD; (*aktu&#xFFFD; (*aktu&#xFFFD; (*aktu&#xFFFD; (*aktu&#xFFFD; (*aktu&#xFFFD; (*aktu&#xFFFD; (*aktu&#xFFFD; (*aktu&#xFFFD; (*aktu&#xFFFD; (*aktu&#xFFFD; (*aktu&#xFFFD; (*aktu&#xFFFD; (*aktu&#xFFFD; (*aktu&#xFFFD; (*aktu&#xFFFD; (*aktu&#xFFFD; (*aktu&#xFFFD; (*aktu&#xFFFD; (*aktu&#xFFFD; (*aktu&#xFFFD; (*aktu&#xFFFD; (*aktu&#xFFFD; (*aktu&#xFFFD; (*aktu&#xFFFD; (*aktu&#xFFFD; (*aktu&#xFFFD; (*aktu&#xFFFD; (*aktu&#xFFFD; (*aktu&#xFFFD; (*aktu&#xFFFD; (*aktu&#xFFFD; (*aktu&#xFFFD; (*aktu&#xFFFD; (*aktu&#xFFFD; (*aktu&#xFFFD; (*aktu&#xFFFD; (*aktu&#xFFFD; (*aktu&#xFFFD; (*aktu&#xFFFD; (*aktu&#xFFFD; (*aktu&#xFFFD; (*aktu&#xFFFD; (*aktu&#xFFFD; (*aktu&#xFFFD; (*aktu&#xFFFD; (*aktu&#xFFFD; (*aktu&#xFFFD; (*aktu&#xFFFD; (*aktu&#xFFFD; (*aktu&#xFFFD; (*aktu&#xFFFD; (*aktu&#xFFFD; (*aktu&#xFFFD; (*aktu&#xFFFD; (*aktu&#xFFFD; (*aktu&#xFFFD; (*aktu&#xFFFD; (*aktu&#xFFFD; (*aktu&#xFFFD; (*aktu&#xFFFD; (*aktu&#xFFFD; (*aktu&#xFFFD; (*aktu&#xFFFD; (*aktu&#xFFFD; (*aktu&#xFFFD; (*aktu&#xFFFD; (*aktu&#xFFFD; (*aktu&#xFFFD; (*aktu&#xFFFD; (*aktu&#xFFFD; (*aktu&#xFFFD; (*aktu&#xFFFD; (*aktu&#xFFFD; (*aktu&#xFFFD; (*aktu&#xFFFD; (*aktu&#xFFFD; (*aktu&#xFFFD; (*aktu&#xFFFD; (*aktu&#xFFFD; (*aktu&#xFFFD; (*aktu&#xFFFD; (*aktu&#xFFFD; (*aktu&#xFFFD; (*aktu&#xFFFD; (*aktu&#xFFFD; (*aktu&#xFFFD; (*aktu&#xFFFD; (*aktu&#xFFFD; (*aktu&#xFFFD; (*aktu&#xFFFD; (*aktu&#xFFFD; (*aktu&#xFFFD; (*aktu&#xFFFD; (*aktu&#xFFFD; (*aktu&#xFFFD; (*aktu&#xFFFD; (*aktu&#xFFFD; (*aktu&#xFFFD; (*aktu&#xFFFD; (*aktu&#xFFFD; (*aktu&#xFFFD; (*aktu&#xFFFD; (*aktu&#xFFFD; (*aktu&#xFFFD; (*aktu&#xFFFD; (*aktu&#xFFFD; (*aktu&#xFFFD; (*aktu&#xFFFD; (*aktu&#xFFFD; (*aktu&#xFFFD; (*aktu&#xFFFD; (*aktu&#xFFFD; (*aktu&#xFFFD; (*aktu&#xFFFD; (*aktu&#xFFFD; (*aktu&#xFFFD; (*aktu&#xFFFD; (*aktu&#xFFFD; (*aktu&#xFFFD; (*aktu&#xFFFD; (*aktu&#xFFFD; (*aktu&#xFFFD; (*aktu&#xFFFD; (*aktu&#xFFFD; (*aktu&#xFFFD; (*aktu&#xFFFD; (*aktu&#xFFFD; (*aktu&#xFFFD; (*aktu&#xFFFD; (*aktu&#xFFFD; (*aktu&#xFFFD; (*aktu&#xFFFD; (*aktu&#xFFFD; (*aktu&#xFFFD; (*aktu&#xFFFD; (*aktu&#xFFFD; (*aktu&#xFFFD; (*aktu&#xFFFD; (*aktu&#xFFFD; (*aktu&#xFFFD; (*aktu&#xFFFD; (*aktu&#xFFFD; (*aktu&#xFFFD; (*aktu&#xFFFD; (*aktu&#xFFFD; (*aktu&#xFFFD; (*aktu&#xFFFD; (*aktu&#xFFFD; (*aktu&#xFFFD; (*aktu&#xFFFD; (*aktu&#xFFFD; (*aktu&#xFFFD; (*aktu&#xFFFD; (*aktu&#xFFFD; (*aktu&#xFFFD; (*aktu&#xFFFD; (*aktu&#xFFFD; (*aktu&#xFFFD; (*aktu&#xFFFD; (*aktu&#xFFFD; (*aktu&#xFFFD; (*aktu&#xFFFD; (*aktu&#xFFFD; (*aktu&#xFFFD; (*aktu&#xFFFD; (*aktu&#xFFFD; (*aktu&#xFFFD; (*aktu&#xFFFD; (*aktu&#xFFFD; (*aktu&#xFFFD; (*aktu&#xFFFD; (*aktu&#xFFFD; (*aktu&#xFFFD; (*aktu&#xFFFD; (*aktu&#xFFFD; (*aktu&#xFFFD; (*aktu&#xFFFD; (*aktu&#xFFFD; (*aktu&#xFFFD; (*aktu&#xFFFD; (*aktu&#xFFFD; (*aktu&#xFFFD; (*aktu&#xFFFD; (*aktu&#xFFFD; (*aktu&#xFFFD; (*aktu&#xFFFD; (*aktu&#xFFFD; (*aktu&#xFFFD; (*aktu&#xFFFD; (*aktu&#xFFFD; (*aktu&#xFFFD; (*aktu&#xFFFD; (*aktu&#xFFFD; (*aktu&#xFFFD; (*aktu&#xFFFD; (*aktu&#xFFFD; (*aktu&#xFFFD; (*aktu&#xFFFD; (*aktu&#xFFFD; (*aktu&#xFFFD; (*aktu&#xFFFD; (*aktu&#xFFFD; (*aktu&#xFFFD; (*aktu&#xFFFD; (*aktu&#xFFFD; (*aktu&#xFFFD; (*aktu&#xFFFD; (*aktu&#xFFFD; (*aktu&#xFFFD; (*aktu&#xFFFD; (*aktu&#xFFFD; (*aktu&#xFFFD; (*aktu&#xFFFD; (*aktu&#xFFFD; (*aktu&#xFFFD; (*aktu&#xFFFD; (*aktu&#xFFFD; (*aktu&#xFFFD; (*aktu&#xFFFD; (*aktu&#xFFFD; (*aktu&#xFFFD; (*aktu&#xFFFD; (*aktu&#xFFFD; (*aktu&#xFFFD; (*aktu&#xFFFD; (*aktu&#xFFFD; (*aktu&#xFFFD; (*aktu&#xFFFD; (*aktu&#xFFFD; (*aktu&#xFFFD; (*aktu&#xFFFD; (*aktu&#xFFFD; (*aktu&#xFFFD; (*aktu&#xFFFD; (*aktu&#xFFFD; (*aktu&#xFFFD; (*aktu&#xFFFD; (*aktu&#xFFFD; (*aktu&#xFFFD; (*aktu&#xFFFD; (*aktu&#xFFFD; (*aktu&#xFFFD; (*aktu&#xFFFD; (*aktu&#xFFFD; (*aktu&#xFFFD; (*aktu&#xFFFD; (*aktu&#xFFFD; (*aktu&#xFFFD; (*aktu&#xFFFD; (*aktu&#xFFFD; (*aktu&#xFFFD; (*aktu&#xFFFD; (*aktu&#xFFFD; (*aktu&#xFFFD; (*aktu&#xFFFD; (*aktu&#xFFFD; (*aktu&#xFFFD; (*aktu&#xFFFD; (*aktu&#xFFFD; (*aktu&#xFFFD; (*aktu&#xFFFD; (*aktu&#xFFFD; (*aktu&#xFFFD; (*aktu&#xFFFD; (*aktu&#xFFFD; (*aktu&#xFFFD; (*aktu&#xFFFD; (*aktu&#xFFFD; (*aktu&#xFFFD; (*aktu&#xFFFD; (*aktu&#xFFFD; (*aktu&#xFFFD; (*aktu&#xFFFD; (*aktu&#xFFFD; (*aktu&#xFFFD; (*aktu&#xFFFD; (*aktu&#xFFFD; (*aktu&#xFFFD; (*aktu&#xFFFD; (*aktu&#xFFFD; (*aktu&#xFFFD; (*aktu&#xFFFD; (*aktu&#xFFFD; (*aktu&#xFFFD; (*aktu&#xFFFD; (*aktu&#xFFFD; (*aktu&#xFFFD; (*aktu&#xFFFD; (*aktu&#xFFFD; (*aktu&#xFFFD; (*aktu&#xFFFD; (*aktu&#xFFFD; (*aktu&#xFFFD; (*aktu&#xFFFD; (*aktu&#xFFFD; (*aktu&#xFFFD; (*aktu&#xFFFD; (*aktu&#xFFFD; (*aktu&#xFFFD; (*aktu&#xFFFD; (*aktu&#xFFFD; (*aktu&#xFFFD; (*aktu&#xFFFD; (*aktu&#xFFFD; (*aktu&#xFFFD; (*aktu&#xFFFD; (*aktu&#xFFFD; (*aktu&#xFFFD; (*aktu&#xFFFD; (*aktu&#xFFFD; (*aktu&#xFFFD; (*aktu&#xFFFD; (*aktu&#xFFFD; (*aktu&#xFFFD; (*aktu&#xFFFD; (*aktu&#xFFFD; (*aktu&#xFFFD; (*aktu&#xFFFD; (*aktu&#xFFFD; (*aktu&#xFFFD; (*aktu&#xFFFD; (*aktu&#xFFFD; (*aktu&#xFFFD; (*aktu&#xFFFD; (*aktu&#xFFFD; (*aktu&#xFFFD; (*aktu&#xFFFD; (*aktu&#xFFFD; (*aktu&#xFFFD; (*aktu&#xFFFD; (*aktu&#xFFFD; (*aktu&#xFFFD; (*aktu&#xFFFD; (*aktu&#xFFFD; (*aktu&#xFFFD; (*aktu&#xFFFD; (*aktu&#xFFFD; (*aktu&#xFFFD; (*aktu&#xFFFD; (*aktu&#xFFFD; (*aktu&#xFFFD; (*aktu&#xFFFD; (*aktu&#xFFFD; (*aktu&#xFFFD; (*aktu&#xFFFD; (*aktu&#xFFFD; (*aktu&#xFFFD; (*aktu&#xFFFD; (*aktu&#xFFFD; (*aktu&#xFFFD; (*aktu&#xFFFD; (*aktu&#xFFFD; (*aktu&#xFFFD; (*aktu&#xFFFD; (*aktu&#xFFFD; (*aktu&#xFFFD; (*aktu&#xFFFD; (*aktu&#xFFFD; (*aktu&#xFFFD; (*aktu&#xFFFD; (*aktu&#xFFFD; (*aktu&#xFFFD; (*aktu&#xFFFD; (*aktu&#xFFFD; (*aktu&#xFFFD; (*aktu&#xFFFD; (*aktu&#xFFFD; (*aktu&#xFFFD; (*aktu&#xFFFD; (*aktu&#xFFFD; (*aktu&#xFFFD; (*aktu&#xFFFD; (*aktu&#xFFFD; (*aktu&#xFFFD; (*aktu&#xFFFD; (*aktu&#xFFFD; (*aktu&#xFFFD; (*aktu&#xFFFD; (*aktu&#xFFFD; (*aktu&#xFFFD; (*aktu&#xFFFD; (*aktu&#xFFFD; (*aktu&#xFFFD; (*aktu&#xFFFD; (*aktu&#xFFFD; (*aktu&#xFFFD; (*aktu&#xFFFD; (*aktu&#xFFFD; (*aktu&#xFFFD; (*aktu&#xFFFD; (*aktu&#xFFFD; (*aktu&#xFFFD; (*aktu&#xFFFD; (*aktu&#xFFFD; (*aktu&#xFFFD; (*aktu&#xFFFD; (*aktu&#xFFFD; (*aktu&#xFFFD; (*aktu&#xFFFD; (*aktu&#xFFFD; (*aktu&#xFFFD; (*aktu&#xFFFD; (*aktu&#xFFFD; (*aktu&#xFFFD; (*aktu&#xFFFD; (*aktu&#xFFFD; (*aktu&#xFFFD; (*aktu&#xFFFD; (*aktu&#xFFFD; (*aktu&#xFFFD; (*aktu&#xFFFD; (*aktu&#xFFFD; (*aktu&#xFFFD; (*aktu&#xFFFD; (*aktu&#xFFFD; (*aktu&#xFFFD; (*aktu&#xFFFD; (*aktu&#xFFFD; (*aktu&#xFFFD; (*aktu&#xFFFD; (*aktu&#xFFFD; (*aktu&#xFFFD; (*aktu&#xFFFD; (*aktu&#xFFFD; (*aktu&#xFFFD; (*aktu&#xFFFD; (*aktu&#xFFFD; (*aktu&#xFFFD; (*aktu&#xFFFD; (*aktu&#xFFFD; (*aktu&#xFFFD; (*aktu&#xFFFD; (*aktu&#xFFFD; (*aktu&#xFFFD; (*aktu&#xFFFD; (*aktu&#xFFFD; (*aktu&#xFFFD; (*aktu&#xFFFD; (*aktu&#xFFFD; (*aktu&#xFFFD; (*aktu&#xFFFD; (*aktu&#xFFFD; (*aktu&#xFFFD; (*aktu&#xFFFD; (*aktu&#xFFFD; (*aktu&#xFFFD; (*aktu&#xFFFD; (*aktu&#xFFFD; (*aktu&#xFFFD; (*aktu&#xFFFD; (*aktu&#xFFFD; (*aktu&#xFFFD; (*aktu&#xFFFD; (*aktu&#xFFFD; (*aktu&#xFFFD; (*aktu&#xFFFD; (*aktu&#xFFFD; (*aktu&#xFFFD; (*aktu&#xFFFD; (*aktu&#xFFFD; (*aktu&#xFFFD; (*aktu&#xFFFD; (*aktu&#xFFFD; (*aktu&#xFFFD; (*aktu&#xFFFD; (*aktu&#xFFFD; (*aktu&#xFFFD; (*aktu&#xFFFD; (*aktu&#xFFFD; (*aktu&#xFFFD; (*aktu&#xFFFD; (*aktu&#xFFFD; (*aktu&#xFFFD; (*aktu&#xFFFD; (*aktu&#xFFFD; (*aktu&#xFFFD; (*aktu&#xFFFD; (*aktu&#xFFFD; (*aktu&#xFFFD; (*aktu&#xFFFD; (*aktu&#xFFFD; (*aktu&#xFFFD; (*aktu&#xFFFD; (*aktu&#xFFFD; (*aktu&#xFFFD; (*aktu&#xFFFD; (*aktu&#xFFFD; (*aktu&#xFFFD; (*aktu&#xFFFD; (*aktu&#xFFFD; (*aktu&#xFFFD; (*aktu&#xFFFD; (*aktu&#xFFFD; (*aktu&#xFFFD; (*aktu&#xFFFD; (*aktu&#xFFFD; (*aktu&#xFFFD; (*aktu&#xFFFD; (*aktu&#xFFFD; (*aktu&#xFFFD; (*aktu&#xFFFD; (*aktu&#xFFFD; (*aktu&#xFFFD; (*aktu&#xFFFD; (*aktu&#xFFFD; (*aktu&#xFFFD; (*aktu&#xFFFD; (*aktu&#xFFFD; (*aktu&#xFFFD; (*aktu&#xFFFD; (*aktu&#xFFFD; (*aktu&#xFFFD; (*aktu&#xFFFD; (*aktu&#xFFFD; (*aktu&#xFFFD; (*aktu&#xFFFD; (*aktu&#xFFFD; (*aktu&#xFFFD; (*aktu&#xFFFD; (*aktu&#xFFFD; (*aktu&#xFFFD; (*aktu&#xFFFD; (*aktu&#xFFFD; (*aktu&#xFFFD; (*aktu&#xFFFD; (*aktu&#xFFFD; (*aktu&#xFFFD; (*aktu&#xFFFD; (*aktu&#xFFFD; (*aktu&#xFFFD; (*aktu&#xFFFD; (*aktu&#xFFFD; (*aktu&#xFFFD; (*aktu&#xFFFD; (*aktu&#xFFFD; (*aktu&#xFFFD; (*aktu&#xFFFD; (*aktu&#xFFFD; (*aktu&#xFFFD; (*aktu&#xFFFD; (*aktu&#xFFFD; (*aktu&#xFFFD; (*aktu&#xFFFD; (*aktu&#xFFFD; (*aktu&#xFFFD; (*aktu&#xFFFD; (*aktu&#xFFFD; (*aktu&#xFFFD; (*aktu&#xFFFD; (*aktu&#xFFFD; (*aktu&#xFFFD; (*aktu&#xFFFD; (*aktu&#xFFFD; (*aktu&#xFFFD; (*aktu&#xFFFD; (*aktu&#xFFFD; (*aktu&#xFFFD; (*aktu&#xFFFD; (*aktu&#xFFFD; (*aktu&#xFFFD; (*aktu&#xFFFD; (*aktu&#xFFFD; (*aktu&#xFFFD; (*aktu&#xFFFD; (*aktu&#xFFFD; (*aktu&#xFFFD; (*aktu&#xFFFD; (*aktu&#xFFFD; (*aktu&#xFFFD; (*aktu&#xFFFD; (*aktu&#xFFFD; (*aktu&#xFFFD; (*aktu&#xFFFD; (*aktu&#xFFFD; (*aktu&#xFFFD; (*aktu&#xFFFD; (*aktu&#xFFFD; (*aktu&#xFFFD; (*aktu&#xFFFD; (*aktu&#xFFFD; (*aktu&#xFFFD; (*aktu&#xFFFD; (*aktu&#xFFFD; (*aktu&#xFFFD; (*aktu&#xFFFD; (*aktu&#xFFFD; (*aktu&#xFFFD; (*aktu&#xFFFD; (*aktu&#xFFFD; (*aktu&#xFFFD; (*aktu&#xFFFD; (*aktu&#xFFFD; (*aktu&#xFFFD; (*aktu&#xFFFD; (*aktu&#xFFFD; (*aktu&#xFFFD; (*aktu&#xFFFD; (*aktu&#xFFFD; (*aktu&#xFFFD; (*aktu&#xFFFD; (*aktu&#xFFFD; (*aktu&#xFFFD; (*aktu&#xFFFD; (*aktu&#xFFFD; (*aktu&#xFFFD; (*aktu&#xFFFD; (*aktu&#xFFFD; (*aktu&#xFFFD; (*aktu&#xFFFD; (*aktu&#xFFFD; (*aktu&#xFFFD; (*aktu&#xFFFD; (*aktu&#xFFFD; (*aktu&#xFFFD; (*aktu&#xFFFD; (*aktu&#xFFFD; (*aktu&#xFFFD; (*aktu&#xFFFD; (*aktu&#xFFFD; (*aktu&#xFFFD; (*aktu&#xFFFD; (*aktu&#xFFFD; (*aktu&#xFFFD; (*aktu&#xFFFD; (*aktu&#xFFFD; (*aktu&#xFFFD; (*aktu&#xFFFD; (*aktu&#xFFFD; (*aktu&#xFFFD; (*aktu&#xFFFD; (*aktu&#xFFFD; (*aktu&#xFFFD; (*aktu&#xFFFD; (*aktu&#xFFFD; (*aktu&#xFFFD; (*aktu&#xFFFD; (*aktu&#xFFFD; (*aktu&#xFFFD; (*aktu&#xFFFD; (*aktu&#xFFFD; (*aktu&#xFFFD; (*aktu&#xFFFD; (*aktu&#xFFFD; (*aktu&#xFFFD; (*aktu&#xFFFD; (*aktu&#xFFFD; (*aktu&#xFFFD; (*aktu&#xFFFD; (*aktu&#xFFFD; (*aktu&#xFFFD; (*aktu&#xFFFD; (*aktu&#xFFFD; (*aktu&#xFFFD; (*aktu&#xFFFD; (*aktu&#xFFFD; (*aktu&#xFFFD; (*aktu&#xFFFD; (*aktu&#xFFFD; (*aktu&#xFFFD; (*aktu&#xFFFD; (*aktu&#xFFFD; (*aktu&#xFFFD; (*aktu&#xFFFD; (*aktu&#xFFFD; (*aktu&#xFFFD; (*aktu&#xFFFD; (*aktu&#xFFFD; (*aktu&#xFFFD; (*aktu&#xFFFD; (*aktu&#xFFFD; (*aktu&#xFFFD; (*aktu&#xFFFD; (*aktu&#xFFFD; (*aktu&#xFFFD; (*aktu&#xFFFD; (*aktu&#xFFFD; (*aktu&#xFFFD; (*aktu&#xFFFD; (*aktu&#xFFFD; (*aktu&#xFFFD; (*aktu&#xFFFD; (*aktu&#xFFFD; (*aktu&#xFFFD; (*aktu&#xFFFD; (*aktu&#xFFFD; (*aktu&#xFFFD; (*aktu&#xFFFD; (*aktu&#xFFFD; (*aktu&#xFFFD; (*aktu&#xFFFD; (*aktu&#xFFFD; (*aktu&#xFFFD; (*aktu&#xFFFD; (*aktu&#xFFFD; (*aktu&#xFFFD; (*aktu&#xFFFD; (*aktu&#xFFFD; (*aktu&#xFFFD; (*aktu&#xFFFD; (*aktu&#xFFFD; (*aktu&#xFFFD; (*aktu&#xFFFD; (*aktu&#xFFFD; (*aktu&#xFFFD; (*aktu&#xFFFD; (*aktu&#xFFFD; (*aktu&#xFFFD; (*aktu&#xFFFD; (*aktu&#xFFFD; (*aktu&#xFFFD; (*aktu&#xFFFD; (*aktu&#xFFFD; (*aktu&#xFFFD; (*aktu&#xFFFD; (*aktu&#xFFFD; (*aktu&#xFFFD; (*aktu&#xFFFD; (*aktu&#xFFFD; (*aktu&#xFFFD; (*aktu&#xFFFD; (*aktu&#xFFFD; (*aktu&#xFFFD; (*aktu&#xFFFD; (*aktu&#xFFFD; (*aktu&#xFFFD; (*aktu&#xFFFD; (*aktu&#xFFFD; (*aktu&#xFFFD; (*aktu&#xFFFD; (*aktu&#xFFFD; (*aktu&#xFFFD; (*aktu&#xFFFD; (*aktu&#xFFFD; (*aktu&#xFFFD; (*aktu&#xFFFD; (*aktu&#xFFFD; (*aktu&#xFFFD; (*aktu&#xFFFD; (*aktu&#xFFFD; (*aktu&#xFFFD; (*aktu&#xFFFD; (*aktu&#xFFFD; (*aktu&#xFFFD; (*aktu&#xFFFD; (*aktu&#xFFFD; (*aktu&#xFFFD; (*aktu&#xFFFD; (*aktu&#xFFFD; (*aktu&#xFFFD; (*aktu&#xFFFD; (*aktu&#xFFFD; (*aktu&#xFFFD; (*aktu&#xFFFD; (*aktu&#xFFFD; (*aktu&#xFFFD; (*aktu&#xFFFD; (*aktu&#xFFFD; (*aktu&#xFFFD; (*aktu&#xFFFD; (*aktu&#xFFFD; (*aktu&#xFFFD; (*aktu&#xFFFD; (*aktu&#xFFFD; (*aktu&#xFFFD; (*aktu&#xFFFD; (*aktu&#xFFFD; (*aktu&#xFFFD; (*aktu&#xFFFD; (*aktu&#xFFFD; (*aktu&#xFFFD; (*aktu&#xFFFD; (*aktu&#xFFFD; (*aktu&#xFFFD; (*aktu&#xFFFD; (*aktu&#xFFFD; (*aktu&#xFFFD; (*aktu&#xFFFD; (*aktu&#xFFFD; (*aktu&#xFFFD; (*aktu&#xFFFD; (*aktu&#xFFFD; (*aktu&#xFFFD; (*aktu&#xFFFD; (*aktu&#xFFFD; (*aktu&#xFFFD; (*aktu&#xFFFD; (*aktu&#xFFFD; (*aktu&#xFFFD; (*aktu&#xFFFD; (*aktu&#xFFFD; (*aktu&#xFFFD; (*aktu&#xFFFD; (*aktu&#xFFFD; (*aktu&#xFFFD; (*aktu&#xFFFD; (*aktu&#xFFFD; (*aktu&#xFFFD; (*aktu&#xFFFD; (*aktu&#xFFFD; (*aktu&#xFFFD; (*aktu&#xFFFD; (*aktu&#xFFFD; (*aktu&#xFFFD; (*aktu&#xFFFD; (*aktu&#xFFFD; (*aktu&#xFFFD; (*aktu&#xFFFD; (*aktu&#xFFFD; (*aktu&#xFFFD; (*aktu&#xFFFD; (*aktu&#xFFFD; (*aktu&#xFFFD; (*aktu&#xFFFD; (*aktu&#xFFFD; (*aktu&#xFFFD; (*aktu&#xFFFD; (*aktu&#xFFFD; (*aktu&#xFFFD; (*aktu&#xFFFD; (*aktu&#xFFFD; (*aktu&#xFFFD; (*aktu&#xFFFD; (*aktu&#xFFFD; (*aktu&#xFFFD; (*aktu&#xFFFD; (*aktu&#xFFFD; (*aktu&#xFFFD; (*aktu&#xFFFD; (*aktu&#xFFFD; (*aktu&#xFFFD; (*aktu&#xFFFD; (*aktu&#xFFFD; (*aktu&#xFFFD; (*aktu&#xFFFD; (*aktu&#xFFFD; (*aktu&#xFFFD; (*aktu&#xFFFD; (*aktu&#xFFFD; (*aktu&#xFFFD; (*aktu&#xFFFD; (*aktu&#xFFFD; (*aktu&#xFFFD; (*aktu&#xFFFD; (*aktu&#xFFFD; (*aktu&#xFFFD; (*aktu&#xFFFD; (*aktu&#xFFFD; (*aktu&#xFFFD; (*aktu&#xFFFD; (*aktu&#xFFFD; (*aktu&#xFFFD; (*aktu&#xFFFD; (*aktu&#xFFFD; (*aktu&#xFFFD; (*aktu&#xFFFD; (*aktu&#xFFFD; (*aktu&#xFFFD; (*aktu&#xFFFD; (*aktu&#xFFFD; (*aktu&#xFFFD; (*aktu&#xFFFD; (*aktu&#xFFFD; (*aktu&#xFFFD; (*aktu&#xFFFD; (*aktu&#xFFFD; (*aktu&#xFFFD; (*aktu&#xFFFD; (*aktu&#xFFFD; (*aktu&#xFFFD; (*aktu&#xFFFD; (*aktu&#xFFFD; (*aktu&#xFFFD; (*aktu&#xFFFD; (*aktu&#xFFFD; (*aktu&#xFFFD; (*aktu&#xFFFD; (*aktu&#xFFFD; (*aktu&#xFFFD; (*aktu&#xFFFD; (*aktu&#xFFFD; (*aktu&#xFFFD; (*aktu&#xFFFD; (*aktu&#xFFFD; (*aktu&#xFFFD; (*aktu&#xFFFD; (*aktu&#xFFFD; (*aktu&#xFFFD; (*aktu&#xFFFD; (*aktu&#xFFFD; (*aktu&#xFFFD; (*aktu&#xFFFD; (*aktu&#xFFFD; (*aktu&#xFFFD; (*aktu&#xFFFD; (*aktu&#xFFFD; (*aktu&#xFFFD; (*aktu&#xFFFD; (*aktu&#xFFFD; (*aktu&#xFFFD; (*aktu&#xFFFD; (*aktu&#xFFFD; (*aktu&#xFFFD; (*aktu&#xFFFD; (*aktu&#xFFFD; (*aktu&#xFFFD; (*aktu&#xFFFD; (*aktu&#xFFFD; (*aktu&#xFFFD; (*aktu&#xFFFD; (*aktu&#xFFFD; (*aktu&#xFFFD; (*aktu&#xFFFD; (*aktu&#xFFFD; (*aktu&#xFFFD; (*aktu&#xFFFD; (*aktu&#xFFFD; (*aktu&#xFFFD; (*aktu&#xFFFD; (*aktu&#xFFFD; (*aktu&#xFFFD; (*aktu&#xFFFD; (*aktu&#xFFFD; (*aktu&#xFFFD; (*aktu&#xFFFD; (*aktu&#xFFFD; (*aktu&#xFFFD; (*aktu&#xFFFD; (*aktu&#xFFFD; (*aktu&#xFFFD; (*aktu&#xFFFD; (*aktu&#xFFFD; (*aktu&#xFFFD; (*aktu&#xFFFD; (*aktu&#xFFFD; (*aktu&#xFFFD; (*aktu&#xFFFD; (*aktu&#xFFFD; (*aktu&#xFFFD; (*aktu&#xFFFD; (*aktu&#xFFFD; (*aktu&#xFFFD; (*aktu&#xFFFD; (*aktu&#xFFFD; (*aktu&#xFFFD; (*aktu&#xFFFD; (*aktu&#xFFFD; (*aktu&#xFFFD; (*aktu&#xFFFD; (*aktu&#xFFFD; (*aktu&#xFFFD; (*aktu&#xFFFD; (*aktu&#xFFFD; (*aktu&#xFFFD; (*aktu&#xFFFD; (*aktu&#xFFFD; (*aktu&#xFFFD; (*aktu&#xFFFD; (*aktu&#xFFFD; (*aktu&#xFFFD; (*aktu&#xFFFD; (*aktu&#xFFFD; (*aktu&#xFFFD; (*aktu&#xFFFD; (*aktu&#xFFFD; (*aktu&#xFFFD; (*aktu&#xFFFD; (*aktu&#xFFFD; (*aktu&#xFFFD; (*aktu&#xFFFD; (*aktu&#xFFFD; (*aktu&#xFFFD; (*aktu&#xFFFD; (*aktu&#xFFFD; (*aktu&#xFFFD; (*aktu&#xFFFD; (*aktu&#xFFFD; (*aktu&#xFFFD; (*aktu&#xFFFD; (*aktu&#xFFFD; (*aktu&#xFFFD; (*aktu&#xFFFD; (*aktu&#xFFFD; (*aktu&#xFFFD; (*aktu&#xFFFD; (*aktu&#xFFFD; (*aktu&#xFFFD; (*aktu&#xFFFD; (*aktu&#xFFFD; (*aktu&#xFFFD; (*aktu&#xFFFD; (*aktu&#xFFFD; (*aktu&#xFFFD; (*aktu&#xFFFD; (*aktu&#xFFFD; (*aktu&#xFFFD; (*aktu&#xFFFD; (*aktu&#xFFFD; (*aktu&#xFFFD; (*aktu&#xFFFD; (*aktu&#xFFFD; (*aktu&#xFFFD; (*aktu&#xFFFD; (*aktu&#xFFFD; (*aktu&#xFFFD; (*aktu&#xFFFD; (*aktu&#xFFFD; (*aktu&#xFFFD; (*aktu&#xFFFD; (*aktu&#xFFFD; (*aktu&#xFFFD; (*aktu&#xFFFD; (*aktu&#xFFFD; (*aktu&#xFFFD; (*aktu&#xFFFD; (*aktu&#xFFFD; (*aktu&#xFFFD; (*aktu&#xFFFD; (*aktu&#xFFFD; (*aktu&#xFFFD; (*aktu&#xFFFD; (*aktu&#xFFFD; (*aktu&#xFFFD; (*aktu&#xFFFD; (*aktu&#xFFFD; (*aktu&#xFFFD; (*aktu&#xFFFD; (*aktu&#xFFFD; (*aktu&#xFFFD; (*aktu&#xFFFD; (*aktu&#xFFFD; (*aktu&#xFFFD; (*aktu&#xFFFD; (*aktu&#xFFFD; (*aktu&#xFFFD; (*aktu&#xFFFD; (*aktu&#xFFFD; (*aktu&#xFFFD; (*aktu&#xFFFD; (*aktu&#xFFFD; (*aktu&#xFFFD; (*aktu&#xFFFD; (*aktu&#xFFFD; (*aktu&#xFFFD; (*aktu&#xFFFD; (*aktu&#xFFFD; (*aktu&#xFFFD; (*aktu&#xFFFD; (*aktu&#xFFFD; (*aktu&#xFFFD; (*aktu&#xFFFD; (*aktu&#xFFFD; (*aktu&#xFFFD; (*aktu&#xFFFD; (*aktu&#xFFFD; (*aktu&#xFFFD; (*aktu&#xFFFD; (*aktu&#xFFFD; (*aktu&#xFFFD; (*aktu&#xFFFD; (*aktu&#xFFFD; (*aktu&#xFFFD; (*aktu&#xFFFD; (*aktu&#xFFFD; (*aktu&#xFFFD; (*aktu&#xFFFD; (*aktu&#xFFFD; (*aktu&#xFFFD; (*aktu&#xFFFD; (*aktu&#xFFFD; (*aktu&#xFFFD; (*aktu&#xFFFD; (*aktu&#xFFFD; (*aktu&#xFFFD; (*aktu&#xFFFD; (*aktu&#xFFFD; (*aktu&#xFFFD; (*aktu&#xFFFD; (*aktu&#xFFFD; (*aktu&#xFFFD; (*aktu&#xFFFD; (*aktu&#xFFFD; (*aktu&#xFFFD; (*aktu&#xFFFD; (*aktu&#xFFFD; (*aktu&#xFFFD; (*aktu&#xFFFD; (*aktu&#xFFFD; (*aktu&#xFFFD; (*aktu&#xFFFD; (*aktu&#xFFFD; (*aktu&#xFFFD; (*aktu&#xFFFD; (*aktu&#xFFFD; (*aktu&#xFFFD; (*aktu&#xFFFD; (*aktu&#xFFFD; (*aktu&#xFFFD; (*aktu&#xFFFD; (*aktu&#xFFFD; (*aktu&#xFFFD; (*aktu&#xFFFD; (*aktu&#xFFFD; (*aktu&#xFFFD; (*aktu&#xFFFD; (*aktu&#xFFFD; (*aktu&#xFFFD; (*aktu&#xFFFD; (*aktu&#xFFFD; (*aktu&#xFFFD; (*aktu&#xFFFD; (*aktu&#xFFFD; (*aktu&#xFFFD; (*aktu&#xFFFD; (*aktu&#xFFFD; (*aktu&#xFFFD; (*aktu&#xFFFD; (*aktu&#xFFFD; (*aktu&#xFFFD; (*aktu&#xFFFD; (*aktu&#xFFFD; (*aktu&#xFFFD; (*aktu&#xFFFD; (*aktu&#xFFFD; (*aktu&#xFFFD; (*aktu&#xFFFD; (*aktu&#xFFFD; (*aktu&#xFFFD; (*aktu&#xFFFD; (*aktu&#xFFFD; (*aktu&#xFFFD; (*aktu&#xFFFD; (*aktu&#xFFFD; (*aktu&#xFFFD; (*aktu&#xFFFD; (*aktu&#xFFFD; (*aktu&#xFFFD; (*aktu&#xFFFD; (*aktu&#xFFFD; (*aktu&#xFFFD; (*aktu&#xFFFD; (*aktu&#xFFFD; (*aktu&#xFFFD; (*aktu&#xFFFD; (*aktu&#xFFFD; (*aktu&#xFFFD; (*aktu&#xFFFD; (*aktu&#xFFFD; (*aktu&#xFFFD; (*aktu&#xFFFD; (*aktu&#xFFFD; (*aktu&#xFFFD; (*aktu&#xFFFD; (*aktu&#xFFFD; (*aktu&#xFFFD; (*aktu&#xFFFD; (*aktu&#xFFFD; (*aktu&#xFFFD; (*aktu&#xFFFD; (*aktu&#xFFFD; (*aktu&#xFFFD; (*aktu&#xFFFD; (*aktu&#xFFFD; (*aktu&#xFFFD; (*aktu&#xFFFD; (*aktu&#xFFFD; (*aktu&#xFFFD; (*aktu&#xFFFD; (*aktu&#xFFFD; (*aktu&#xFFFD; (*aktu&#xFFFD; (*aktu&#xFFFD; (*aktu&#xFFFD; (*aktu&#xFFFD; (*aktu&#xFFFD; (*aktu&#xFFFD; (*aktu&#xFFFD; (*aktu&#xFFFD; (*aktu&#xFFFD; (*aktu&#xFFFD; (*aktu&#xFFFD; (*aktu&#xFFFD; (*aktu&#xFFFD; (*aktu&#xFFFD; (*aktu&#xFFFD; (*aktu&#xFFFD; (*aktu&#xFFFD; (*aktu&#xFFFD; (*aktu&#xFFFD; (*aktu&#xFFFD; (*aktu&#xFFFD; (*aktu&#xFFFD; (*aktu&#xFFFD; (*aktu&#xFFFD; (*aktu&#xFFFD; (*aktu&#xFFFD; (*aktu&#xFFFD; (*aktu&#xFFFD; (*aktu&#xFFFD; (*aktu&#xFFFD; (*aktu&#xFFFD; (*aktu&#xFFFD; (*aktu&#xFFFD; (*aktu&#xFFFD; (*aktu&#xFFFD; (*aktu&#xFFFD; (*aktu&#xFFFD; (*aktu&#xFFFD; (*aktu&#xFFFD; (*aktu&#xFFFD; (*aktu&#xFFFD; (*aktu&#xFFFD; (*aktu&#xFFFD; (*aktu&#xFFFD; (*aktu&#xFFFD; (*aktu&#xFFFD; (*aktu&#xFFFD; (*aktu&#xFFFD; (*aktu&#xFFFD; (*aktu&#xFFFD; (*aktu&#xFFFD; (*aktu&#xFFFD; (*aktu&#xFFFD; (*aktu&#xFFFD; (*aktu&#xFFFD; (*aktu&#xFFFD; (*aktu&#xFFFD; (*aktu&#xFFFD; (*aktu&#xFFFD; (*aktu&#xFFFD; (*aktu&#xFFFD; (*aktu&#xFFFD; (*aktu&#xFFFD; (*aktu&#xFFFD; (*aktu&#xFFFD; (*aktu&#xFFFD; (*aktu&#xFFFD; (*aktu&#xFFFD; (*aktu&#xFFFD; (*aktu&#xFFFD; (*aktu&#xFFFD; (*aktu&#xFFFD; (*aktu&#xFFFD; (*aktu&#xFFFD; (*aktu&#xFFFD; (*aktu&#xFFFD; (*aktu&#xFFFD; (*aktu&#xFFFD; (*aktu&#xFFFD; (*aktu&#xFFFD; (*aktu&#xFFFD; (*aktu&#xFFFD; (*aktu&#xFFFD; (*aktu&#xFFFD; (*aktu&#xFFFD; (*aktu&#xFFFD; (*aktu&#xFFFD; (*aktu&#xFFFD; (*aktu&#xFFFD; (*aktu&#xFFFD; (*aktu&#xFFFD; (*aktu&#xFFFD; (*aktu&#xFFFD; (*aktu&#xFFFD; (*aktu&#xFFFD; (*aktu&#xFFFD; (*aktu&#xFFFD; (*aktu&#xFFFD; (*aktu&#xFFFD; (*aktu&#xFFFD; (*aktu&#xFFFD; (*aktu&#xFFFD; (*aktu&#xFFFD; (*aktu&#xFFFD; (*aktu&#xFFFD; (*aktu&#xFFFD; (*aktu&#xFFFD; (*aktu&#xFFFD; (*aktu&#xFFFD; (*aktu&#xFFFD; (*aktu&#xFFFD; (*aktu&#xFFFD; (*aktu&#xFFFD; (*aktu&#xFFFD; (*aktu&#xFFFD; (*aktu&#xFFFD; (*aktu&#xFFFD; (*aktu&#xFFFD; (*aktu&#xFFFD; (*aktu&#xFFFD; (*aktu&#xFFFD; (*aktu&#xFFFD; (*aktu&#xFFFD; (*aktu&#xFFFD; (*aktu&#xFFFD; (*aktu&#xFFFD; (*aktu&#xFFFD; (*aktu&#xFFFD; (*aktu&#xFFFD; (*aktu&#xFFFD; (*aktu&#xFFFD; (*aktu&#xFFFD; (*aktu&#xFFFD; (*aktu&#xFFFD; (*aktu&#xFFFD; (*aktu&#xFFFD; (*aktu&#xFFFD; (*aktu&#xFFFD; (*aktu&#xFFFD; (*aktu&#xFFFD; (*aktu&#xFFFD; (*aktu&#xFFFD; (*aktu&#xFFFD; (*aktu&#xFFFD; (*aktu&#xFFFD; (*aktu&#xFFFD; (*aktu&#xFFFD; (*aktu&#xFFFD; (*aktu&#xFFFD; (*aktu&#xFFFD; (*aktu&#xFFFD; (*aktu&#xFFFD; (*aktu&#xFFFD; (*aktu&#xFFFD; (*aktu&#xFFFD; (*aktu&#xFFFD; (*aktu&#xFFFD; (*aktu&#xFFFD; (*aktu&#xFFFD; (*aktu&#xFFFD; (*aktu&#xFFFD; (*aktu&#xFFFD; (*aktu&#xFFFD; (*aktu&#xFFFD; (*aktu&#xFFFD; (*aktu&#xFFFD; (*aktu&#xFFFD; (*aktu&#xFFFD; (*aktu&#xFFFD; (*aktu&#xFFFD; (*aktu&#xFFFD; (*aktu&#xFFFD; (*aktu&#xFFFD; (*aktu&#xFFFD; (*aktu&#xFFFD; (*aktu&#xFFFD; (*aktu&#xFFFD; (*aktu&#xFFFD; (*aktu&#xFFFD; (*aktu&#xFFFD; (*aktu&#xFFFD; (*aktu&#xFFFD; (*aktu&#xFFFD; (*aktu&#xFFFD; (*aktu&#xFFFD; (*aktu&#xFFFD; (*aktu&#xFFFD; (*aktu&#xFFFD; (*aktu&#xFFFD; (*aktu&#xFFFD; (*aktu&#xFFFD; (*aktu&#xFFFD; (*aktu&#xFFFD; (*aktu&#xFFFD; (*aktu&#xFFFD; (*aktu&#xFFFD; (*aktu&#xFFFD; (*aktu&#xFFFD; (*aktu&#xFFFD; (*aktu&#xFFFD; (*aktu&#xFFFD; (*aktu&#xFFFD; (*aktu&#xFFFD; (*aktu&#xFFFD; (*aktu&#xFFFD; (*aktu&#xFFFD; (*aktu&#xFFFD; (*aktu&#xFFFD; (*aktu&#xFFFD; (*aktu&#xFFFD; (*aktu&#xFFFD; (*aktu&#xFFFD; (*aktu&#xFFFD; (*aktu&#xFFFD; (*aktu&#xFFFD; (*aktu&#xFFFD; (*aktu&#xFFFD; (*aktu&#xFFFD; (*aktu&#xFFFD; (*aktu&#xFFFD; (*aktu&#xFFFD; (*aktu&#xFFFD; (*aktu&#xFFFD; (*aktu&#xFFFD; (*aktu&#xFFFD; (*aktu&#xFFFD; (*aktu&#xFFFD; (*aktu&#xFFFD; (*aktu&#xFFFD; (*aktu&#xFFFD; (*aktu&#xFFFD; (*aktu&#xFFFD; (*aktu&#xFFFD; (*aktu&#xFFFD; (*aktu&#xFFFD; (*aktu&#xFFFD; (*aktu&#xFFFD; (*aktu&#xFFFD; (*aktu&#xFFFD; (*aktu&#xFFFD; (*aktu&#xFFFD; (*aktu&#xFFFD; (*aktu&#xFFFD; (*aktu&#xFFFD; (*aktu&#xFFFD; (*aktu&#xFFFD; (*aktu&#xFFFD; (*aktu&#xFFFD; (*aktu&#xFFFD; (*aktu&#xFFFD; (*aktu&#xFFFD; (*aktu&#xFFFD; (*aktu&#xFFFD; (*aktu&#xFFFD; (*aktu&#xFFFD; (*aktu&#xFFFD; (*aktu&#xFFFD; (*aktu&#xFFFD; (*aktu&#xFFFD; (*aktu&#xFFFD; (*aktu&#xFFFD; (*aktu&#xFFFD; (*aktu&#xFFFD; (*aktu&#xFFFD; (*aktu&#xFFFD; (*aktu&#xFFFD; (*aktu&#xFFFD; (*aktu&#xFFFD; (*aktu&#xFFFD; (*aktu&#xFFFD; (*aktu&#xFFFD; (*aktu&#xFFFD; (*aktu&#xFFFD; (*aktu&#xFFFD; (*aktu&#xFFFD; (*aktu&#xFFFD; (*aktu&#xFFFD; (*aktu&#xFFFD; (*aktu&#xFFFD; (*aktu&#xFFFD; (*aktu&#xFFFD; (*aktu&#xFFFD; (*aktu&#xFFFD; (*aktu&#xFFFD; (*aktu&#xFFFD; (*aktu&#xFFFD; (*aktu&#xFFFD; (*aktu&#xFFFD; (*aktu&#xFFFD; (*aktu&#xFFFD; (*aktu&#xFFFD; (*aktu&#xFFFD; (*aktu&#xFFFD; (*aktu&#xFFFD; (*aktu&#xFFFD; (*aktu&#xFFFD; (*aktu&#xFFFD; (*aktu&#xFFFD; (*aktu&#xFFFD; (*aktu&#xFFFD; (*aktu&#xFFFD; (*aktu&#xFFFD; (*aktu&#xFFFD; (*aktu&#xFFFD; (*aktu&#xFFFD; (*aktu&#xFFFD; (*aktu&#xFFFD; (*aktu&#xFFFD; (*aktu&#xFFFD; (*aktu&#xFFFD; (*aktu&#xFFFD; (*aktu&#xFFFD; (*aktu&#xFFFD; (*aktu&#xFFFD; (*aktu&#xFFFD; (*aktu&#xFFFD; (*aktu&#xFFFD; (*aktu&#xFFFD; (*aktu&#xFFFD; (*aktu&#xFFFD; (*aktu&#xFFFD; (*aktu&#xFFFD; (*aktu&#xFFFD; (*aktu&#xFFFD; (*aktu&#xFFFD; (*aktu&#xFFFD; (*aktu&#xFFFD; (*aktu&#xFFFD; (*aktu&#xFFFD; (*aktu&#xFFFD; (*aktu&#xFFFD; (*aktu&#xFFFD; (*aktu&#xFFFD; (*aktu&#xFFFD; (*aktu&#xFFFD; (*aktu&#xFFFD; (*aktu&#xFFFD; (*aktu&#xFFFD; (*aktu&#xFFFD; (*aktu&#xFFFD; (*aktu&#xFFFD; (*aktu&#xFFFD; (*aktu&#xFFFD; (*aktu&#xFFFD; (*aktu&#xFFFD; (*aktu&#xFFFD; (*aktu&#xFFFD; (*aktu&#xFFFD; (*aktu&#xFFFD; (*aktu&#xFFFD; (*aktu&#xFFFD; (*aktu&#xFFFD; (*aktu&#xFFFD; (*aktu&#xFFFD; (*aktu&#xFFFD; (*aktu&#xFFFD; (*aktu&#xFFFD; (*aktu&#xFFFD; (*aktu&#xFFFD; (*aktu&#xFFFD; (*aktu&#xFFFD; (*aktu&#xFFFD; (*aktu&#xFFFD; (*aktu&#xFFFD; (*aktu&#xFFFD; (*aktu&#xFFFD; (*aktu&#xFFFD; (*aktu&#xFFFD; (*aktu&#xFFFD; (*aktu&#xFFFD; (*aktu&#xFFFD; (*aktu&#xFFFD; (*aktu&#xFFFD; (*aktu&#xFFFD; (*aktu&#xFFFD; (*aktu&#xFFFD; (*aktu&#xFFFD; (*aktu&#xFFFD; (*aktu&#xFFFD; (*aktu&#xFFFD; (*aktu&#xFFFD; (*aktu&#xFFFD; (*aktu&#xFFFD; (*aktu&#xFFFD; (*aktu&#xFFFD; (*aktu&#xFFFD; (*aktu&#xFFFD; (*aktu&#xFFFD; (*aktu&#xFFFD; (*aktu&#xFFFD; (*aktu&#xFFFD; (*aktu&#xFFFD; (*aktu&#xFFFD; (*aktu&#xFFFD; (*aktu&#xFFFD; (*aktu&#xFFFD; (*aktu&#xFFFD; (*aktu&#xFFFD; (*aktu&#xFFFD; (*aktu&#xFFFD; (*aktu&#xFFFD; (*aktu&#xFFFD; (*aktu&#xFFFD; (*aktu&#xFFFD; (*aktu&#xFFFD; (*aktu&#xFFFD; (*aktu&#xFFFD; (*aktu&#xFFFD; (*aktu&#xFFFD; (*aktu&#xFFFD; (*aktu&#xFFFD; (*aktu&#xFFFD; (*aktu&#xFFFD; (*aktu&#xFFFD; (*aktu&#xFFFD; (*aktu&#xFFFD; (*aktu&#xFFFD; (*aktu&#xFFFD; (*aktu&#xFFFD; (*aktu&#xFFFD; (*aktu&#xFFFD; (*aktu&#xFFFD; (*aktu&#xFFFD; (*aktu&#xFFFD; (*aktu&#xFFFD; (*aktu&#xFFFD; (*aktu&#xFFFD; (*aktu&#xFFFD; (*aktu&#xFFFD; (*aktu&#xFFFD; (*aktu&#xFFFD; (*aktu&#xFFFD; (*aktu&#xFFFD; (*aktu&#xFFFD; (*aktu&#xFFFD; (*aktu&#xFFFD; (*aktu&#xFFFD; (*aktu&#xFFFD; (*aktu&#xFFFD; (*aktu&#xFFFD; (*aktu&#xFFFD; (*aktu&#xFFFD; (*aktu&#xFFFD; (*aktu&#xFFFD; (*aktu&#xFFFD; (*aktu&#xFFFD; (*aktu&#xFFFD; (*aktu&#xFFFD; (*aktu&#xFFFD; (*aktu&#xFFFD; (*aktu&#xFFFD; (*aktu&#xFFFD; (*aktu&#xFFFD; (*aktu&#xFFFD; (*aktu&#xFFFD; (*aktu&#xFFFD; (*aktu&#xFFFD; (*aktu&#xFFFD; (*aktu&#xFFFD; (*aktu&#xFFFD; (*aktu&#xFFFD; (*aktu&#xFFFD; (*aktu&#xFFFD; (*aktu&#xFFFD; (*aktu&#xFFFD; (*aktu&#xFFFD; (*aktu&#xFFFD; (*aktu&#xFFFD; (*aktu&#xFFFD; (*aktu&#xFFFD; (*aktu&#xFFFD; (*aktu&#xFFFD; (*aktu&#xFFFD; (*aktu&#xFFFD; (*aktu&#xFFFD; (*aktu&#xFFFD; (*aktu&#xFFFD; (*aktu&#xFFFD; (*aktu&#xFFFD; (*aktu&#xFFFD; (*aktu&#xFFFD; (*aktu&#xFFFD; (*aktu&#xFFFD; (*aktu&#xFFFD; (*aktu&#xFFFD; (*aktu&#xFFFD; (*aktu&#xFFFD; (*aktu&#xFFFD; (*aktu&#xFFFD; (*aktu&#xFFFD; (*aktu&#xFFFD; (*aktu&#xFFFD; (*aktu&#xFFFD; (*aktu&#xFFFD; (*aktu&#xFFFD; (*aktu&#xFFFD; (*aktu&#xFFFD; (*aktu&#xFFFD; (*aktu&#xFFFD; (*aktu&#xFFFD; (*aktu&#xFFFD; (*aktu&#xFFFD; (*aktu&#xFFFD; (*aktu&#xFFFD; (*aktu&#xFFFD; (*aktu&#xFFFD; (*aktu&#xFFFD; (*aktu&#xFFFD; (*aktu&#xFFFD; (*aktu&#xFFFD; (*aktu&#xFFFD; (*aktu&#xFFFD; (*aktu&#xFFFD; (*aktu&#xFFFD; (*aktu&#xFFFD; (*aktu&#xFFFD; (*aktu&#xFFFD; (*aktu&#xFFFD; (*aktu&#xFFFD; (*aktu&#xFFFD; (*aktu&#xFFFD; (*aktu&#xFFFD; (*aktu&#xFFFD; (*aktu&#xFFFD; (*aktu&#xFFFD; (*aktu&#xFFFD; (*aktu&#xFFFD; (*aktu&#xFFFD; (*aktu&#xFFFD; (*aktu&#xFFFD; (*aktu&#xFFFD; (*aktu&#xFFFD; (*aktu&#xFFFD; (*aktu&#xFFFD; (*aktu&#xFFFD; (*aktu&#xFFFD; (*aktu&#xFFFD; (*aktu&#xFFFD; (*aktu&#xFFFD; (*aktu&#xFFFD; (*aktu&#xFFFD; (*aktu&#xFFFD; (*aktu&#xFFFD; (*aktu&#xFFFD; (*aktu&#xFFFD; (*aktu&#xFFFD; (*aktu&#xFFFD; (*aktu&#xFFFD; (*aktu&#xFFFD; (*aktu&#xFFFD; (*aktu&#xFFFD; (*aktu&#xFFFD; (*aktu&#xFFFD; (*aktu&#xFFFD; (*aktu&#xFFFD; (*aktu&#xFFFD; (*aktu&#xFFFD; (*aktu&#xFFFD; (*aktu&#xFFFD; (*aktu&#xFFFD; (*aktu&#xFFFD; (*aktu&#xFFFD; (*aktu&#xFFFD; (*aktu&#xFFFD; (*aktu&#xFFFD; (*aktu&#xFFFD; (*aktu&#xFFFD; (*aktu&#xFFFD; (*aktu&#xFFFD; (*aktu&#xFFFD; (*aktu&#xFFFD; (*aktu&#xFFFD; (*aktu&#xFFFD; (*aktu&#xFFFD; (*aktu&#xFFFD; (*aktu&#xFFFD; (*aktu&#xFFFD; (*aktu&#xFFFD; (*aktu&#xFFFD; (*aktu&#xFFFD; (*aktu&#xFFFD; (*aktu&#xFFFD; (*aktu&#xFFFD; (*aktu&#xFFFD; (*aktu&#xFFFD; (*aktu&#xFFFD; (*aktu&#xFFFD; (*aktu&#xFFFD; (*aktu&#xFFFD; (*aktu&#xFFFD; (*aktu&#xFFFD; (*aktu&#xFFFD; (*aktu&#xFFFD; (*aktu&#xFFFD; (*aktu&#xFFFD; (*aktu&#xFFFD; (*aktu&#xFFFD; (*aktu&#xFFFD; (*aktu&#xFFFD; (*aktu&#xFFFD; (*aktu&#xFFFD; (*aktu&#xFFFD; (*aktu&#xFFFD; (*aktu&#xFFFD; (*aktu&#xFFFD; (*aktu&#xFFFD; (*aktu&#xFFFD; (*aktu&#xFFFD; (*aktu&#xFFFD; (*aktu&#xFFFD; (*aktu&#xFFFD; (*aktu&#xFFFD; (*aktu&#xFFFD; (*aktu&#xFFFD; (*aktu&#xFFFD; (*aktu&#xFFFD; (*aktu&#xFFFD; (*aktu&#xFFFD; (*aktu&#xFFFD; (*aktu&#xFFFD; (*aktu&#xFFFD; (*aktu&#xFFFD; (*aktu&#xFFFD; (*aktu&#xFFFD; (*aktu&#xFFFD; (*aktu&#xFFFD; (*aktu&#xFFFD; (*aktu&#xFFFD; (*aktu&#xFFFD; (*aktu&#xFFFD; (*aktu&#xFFFD; (*aktu&#xFFFD; (*aktu&#xFFFD; (*aktu&#xFFFD; (*aktu&#xFFFD; (*aktu&#xFFFD; (*aktu&#xFFFD; (*aktu&#xFFFD; (*aktu&#xFFFD; (*aktu&#xFFFD; (*aktu&#xFFFD; (*aktu&#xFFFD; (*aktu&#xFFFD; (*aktu&#xFFFD; (*aktu&#xFFFD; (*aktu&#xFFFD; (*aktu&#xFFFD; (*aktu&#xFFFD; (*aktu&#xFFFD; (*aktu&#xFFFD; (*aktu&#xFFFD; (*aktu&#xFFFD; (*aktu&#xFFFD; (*aktu&#xFFFD; (*aktu&#xFFFD; (*aktu&#xFFFD; (*aktu&#xFFFD; (*aktu&#xFFFD; (*aktu&#xFFFD; (*aktu&#xFFFD; (*aktu&#xFFFD; (*aktu&#xFFFD; (*aktu&#xFFFD; (*aktu&#xFFFD; (*aktu&#xFFFD; (*aktu&#xFFFD; (*aktu&#xFFFD; (*aktu&#xFFFD; (*aktu&#xFFFD; (*aktu&#xFFFD; (*aktu&#xFFFD; (*aktu&#xFFFD; (*aktu&#xFFFD; (*aktu&#xFFFD; (*aktu&#xFFFD; (*aktu&#xFFFD; (*aktu&#xFFFD; (*aktu&#xFFFD; (*aktu&#xFFFD; (*aktu&#xFFFD; (*aktu&#xFFFD; (*aktu&#xFFFD; (*aktu&#xFFFD; (*aktu&#xFFFD; (*aktu&#xFFFD; (*aktu&#xFFFD; (*aktu&#xFFFD; (*aktu&#xFFFD; (*aktu&#xFFFD; (*aktu&#xFFFD; (*aktu&#xFFFD; (*aktu&#xFFFD; (*aktu&#xFFFD; (*aktu&#xFFFD; (*aktu&#xFFFD; (*aktu&#xFFFD; (*aktu&#xFFFD; (*aktu&#xFFFD; (*aktu&#xFFFD; (*aktu&#xFFFD; (*aktu&#xFFFD; (*aktu&#xFFFD; (*aktu&#xFFFD; (*aktu&#xFFFD; (*aktu&#xFFFD; (*aktu&#xFFFD; (*aktu&#xFFFD; (*aktu&#xFFFD; (*aktu&#xFFFD; (*aktu&#xFFFD; (*aktu&#xFFFD; (*aktu&#xFFFD; (*aktu&#xFFFD; (*aktu&#xFFFD; (*aktu&#xFFFD; (*aktu&#xFFFD; (*aktu&#xFFFD; (*aktu&#xFFFD; (*aktu&#xFFFD; (*aktu&#xFFFD; (*aktu&#xFFFD; (*aktu&#xFFFD; (*aktu&#xFFFD; (*aktu&#xFFFD; (*aktu&#xFFFD; (*aktu&#xFFFD; (*aktu&#xFFFD; (*aktu&#xFFFD; (*aktu&#xFFFD; (*aktu&#xFFFD; (*aktu&#xFFFD; (*aktu&#xFFFD; (*aktu&#xFFFD; (*aktu&#xFFFD; (*aktu&#xFFFD; (*aktu&#xFFFD; (*aktu&#xFFFD; (*aktu&#xFFFD; (*aktu&#xFFFD; (*aktu&#xFFFD; (*aktu&#xFFFD; (*aktu&#xFFFD; (*aktu&#xFFFD; (*aktu&#xFFFD; (*aktu&#xFFFD; (*aktu&#xFFFD; (*aktu&#xFFFD; (*aktu&#xFFFD; (*aktu&#xFFFD; (*aktu&#xFFFD; (*aktu&#xFFFD; (*aktu&#xFFFD; (*aktu&#xFFFD; (*aktu&#xFFFD; (*aktu&#xFFFD; (*aktu&#xFFFD; (*aktu&#xFFFD; (*aktu&#xFFFD; (*aktu&#xFFFD; (*aktu&#xFFFD; (*aktu&#xFFFD; (*aktu&#xFFFD; (*aktu&#xFFFD; (*aktu&#xFFFD; (*aktu&#xFFFD; (*aktu&#xFFFD; (*aktu&#xFFFD; (*aktu&#xFFFD; (*aktu&#xFFFD; (*aktu&#xFFFD; (*aktu&#xFFFD; (*aktu&#xFFFD; (*aktu&#xFFFD; (*aktu&#xFFFD; (*aktu&#xFFFD; (*aktu&#xFFFD; (*aktu&#xFFFD; (*aktu&#xFFFD; (*aktu&#xFFFD; (*aktu&#xFFFD; (*aktu&#xFFFD; (*aktu&#xFFFD; (*aktu&#xFFFD; (*aktu&#xFFFD; (*aktu&#xFFFD; (*aktu&#xFFFD; (*aktu&#xFFFD; (*aktu&#xFFFD; (*aktu&#xFFFD; (*aktu&#xFFFD; (*aktu&#xFFFD; (*aktu&#xFFFD; (*aktu&#xFFFD; (*aktu&#xFFFD; (*aktu&#xFFFD; (*aktu&#xFFFD; (*aktu&#xFFFD; (*aktu&#xFFFD; (*aktu&#xFFFD; (*aktu&#xFFFD; (*aktu&#xFFFD; (*aktu&#xFFFD; (*aktu&#xFFFD; (*aktu&#xFFFD; (*aktu&#xFFFD; (*aktu&#xFFFD; (*aktu&#xFFFD; (*aktu&#xFFFD; (*aktu&#xFFFD; (*aktu&#xFFFD; (*aktu&#xFFFD; (*aktu&#xFFFD; (*aktu&#xFFFD; (*aktu&#xFFFD; (*aktu&#xFFFD; (*aktu&#xFFFD; (*aktu&#xFFFD; (*aktu&#xFFFD; (*aktu&#xFFFD; (*aktu&#xFFFD; (*aktu&#xFFFD; (*aktu&#xFFFD; (*aktu&#xFFFD; (*aktu&#xFFFD; (*aktu&#xFFFD; (*aktu&#xFFFD; (*aktu&#xFFFD; (*aktu&#xFFFD; (*aktu&#xFFFD; (*aktu&#xFFFD; (*aktu&#xFFFD; (*aktu&#xFFFD; (*aktu&#xFFFD; (*aktu&#xFFFD; (*aktu&#xFFFD; (*aktu&#xFFFD; (*aktu&#xFFFD; (*aktu&#xFFFD; (*aktu&#xFFFD; (*aktu&#xFFFD; (*aktu&#xFFFD; (*aktu&#xFFFD; (*aktu&#xFFFD; (*aktu&#xFFFD; (*aktu&#xFFFD; (*aktu&#xFFFD; (*aktu&#xFFFD; (*aktu&#xFFFD; (*aktu&#xFFFD; (*aktu&#xFFFD; (*aktu&#xFFFD; (*aktu&#xFFFD; (*aktu&#xFFFD; (*aktu&#xFFFD; (*aktu&#xFFFD; (*aktu&#xFFFD; (*aktu&#xFFFD; (*aktu&#xFFFD; (*aktu&#xFFFD; (*aktu&#xFFFD; (*aktu&#xFFFD; (*aktu&#xFFFD; (*aktu&#xFFFD; (*aktu&#xFFFD; (*aktu&#xFFFD; (*aktu&#xFFFD; (*aktu&#xFFFD; (*aktu&#xFFFD; (*aktu&#xFFFD; (*aktu&#xFFFD; (*aktu&#xFFFD; (*aktu&#xFFFD; (*aktu&#xFFFD; (*aktu&#xFFFD; (*aktu&#xFFFD; (*aktu&#xFFFD; (*aktu&#xFFFD; (*aktu&#xFFFD; (*aktu&#xFFFD; (*aktu&#xFFFD; (*aktu&#xFFFD; (*aktu&#xFFFD; (*aktu&#xFFFD; (*aktu&#xFFFD; (*aktu&#xFFFD; (*aktu&#xFFFD; (*aktu&#xFFFD; (*aktu&#xFFFD; (*aktu&#xFFFD; (*aktu&#xFFFD; (*aktu&#xFFFD; (*aktu&#xFFFD; (*aktu&#xFFFD; (*aktu&#xFFFD; (*aktu&#xFFFD; (*aktu&#xFFFD; (*aktu&#xFFFD; (*aktu&#xFFFD; (*aktu&#xFFFD; (*aktu&#xFFFD; (*aktu&#xFFFD; (*aktu&#xFFFD; (*aktu&#xFFFD; (*aktu&#xFFFD; (*aktu&#xFFFD; (*aktu&#xFFFD; (*aktu&#xFFFD; (*aktu&#xFFFD; (*aktu&#xFFFD; (*aktu&#xFFFD; (*aktu&#xFFFD; (*aktu&#xFFFD; (*aktu&#xFFFD; (*aktu&#xFFFD; (*aktu&#xFFFD; (*aktu&#xFFFD; (*aktu&#xFFFD; (*aktu&#xFFFD; (*aktu&#xFFFD; (*aktu&#xFFFD; (*aktu&#xFFFD; (*aktu&#xFFFD; (*aktu&#xFFFD; (*aktu&#xFFFD; (*aktu&#xFFFD; (*aktu&#xFFFD; (*aktu&#xFFFD; (*aktu&#xFFFD; (*aktu&#xFFFD; (*aktu&#xFFFD; (*aktu&#xFFFD; (*aktu&#xFFFD; (*aktu&#xFFFD; (*aktu&#xFFFD; (*aktu&#xFFFD; (*aktu&#xFFFD; (*aktu&#xFFFD; (*aktu&#xFFFD; (*aktu&#xFFFD; (*aktu&#xFFFD; (*aktu&#xFFFD; (*aktu&#xFFFD; (*aktu&#xFFFD; (*aktu&#xFFFD; (*aktu&#xFFFD; (*aktu&#xFFFD; (*aktu&#xFFFD; (*aktu&#xFFFD; (*aktu&#xFFFD; (*aktu&#xFFFD; (*aktu&#xFFFD; (*aktu&#xFFFD; (*aktu&#xFFFD; (*aktu&#xFFFD; (*aktu&#xFFFD; (*aktu&#xFFFD; (*aktu&#xFFFD; (*aktu&#xFFFD; (*aktu&#xFFFD; (*aktu&#xFFFD; (*aktu&#xFFFD; (*aktu&#xFFFD; (*aktu&#xFFFD; (*aktu&#xFFFD; (*aktu&#xFFFD; (*aktu&#xFFFD; (*aktu&#xFFFD; (*aktu&#xFFFD; (*aktu&#xFFFD; (*aktu&#xFFFD; (*aktu&#xFFFD; (*aktu&#xFFFD; (*aktu&#xFFFD; (*aktu&#xFFFD; (*aktu&#xFFFD; (*aktu&#xFFFD; (*aktu&#xFFFD; (*aktu&#xFFFD; (*aktu&#xFFFD; (*aktu&#xFFFD; (*aktu&#xFFFD; (*aktu&#xFFFD; (*aktu&#xFFFD; (*aktu&#xFFFD; (*aktu&#xFFFD; (*aktu&#xFFFD; (*aktu&#xFFFD; (*aktu&#xFFFD; (*aktu&#xFFFD; (*aktu&#xFFFD; (*aktu&#xFFFD; (*aktu&#xFFFD; (*aktu&#xFFFD; (*aktu&#xFFFD; (*aktu&#xFFFD; (*aktu&#xFFFD; (*aktu&#xFFFD; (*aktu&#xFFFD; (*aktu&#xFFFD; (*aktu&#xFFFD; (*aktu&#xFFFD; (*aktu&#xFFFD; (*aktu&#xFFFD; (*aktu&#xFFFD; (*aktu&#xFFFD; (*aktu&#xFFFD; (*aktu&#xFFFD; (*aktu&#xFFFD; (*aktu&#xFFFD; (*aktu&#xFFFD; (*aktu&#xFFFD; (*aktu&#xFFFD; (*aktu&#xFFFD; (*aktu&#xFFFD; (*aktu&#xFFFD; (*aktu&#xFFFD; (*aktu&#xFFFD; (*aktu&#xFFFD; (*aktu&#xFFFD; (*aktu&#xFFFD; (*aktu&#xFFFD; (*aktu&#xFFFD; (*aktu&#xFFFD; (*aktu&#xFFFD; (*aktu&#xFFFD; (*aktu&#xFFFD; (*aktu&#xFFFD; (*aktu&#xFFFD; (*aktu&#xFFFD; (*aktu&#xFFFD; (*aktu&#xFFFD; (*aktu&#xFFFD; (*aktu&#xFFFD; (*aktu&#xFFFD; (*aktu&#xFFFD; (*aktu&#xFFFD; (*aktu&#xFFFD; (*aktu&#xFFFD; (*aktu&#xFFFD; (*aktu&#xFFFD; (*aktu&#xFFFD; (*aktu&#xFFFD; (*aktu&#xFFFD; (*aktu&#xFFFD; (*aktu&#xFFFD; (*aktu&#xFFFD; (*aktu&#xFFFD; (*aktu&#xFFFD; (*aktu&#xFFFD; (*aktu&#xFFFD; (*aktu&#xFFFD; (*aktu&#xFFFD; (*aktu&#xFFFD; (*aktu&#xFFFD; (*aktu&#xFFFD; (*aktu&#xFFFD; (*aktu&#xFFFD; (*aktu&#xFFFD; (*aktu&#xFFFD; (*aktu&#xFFFD; (*aktu&#xFFFD; (*aktu&#xFFFD; (*aktu&#xFFFD; (*aktu&#xFFFD; (*aktu&#xFFFD; (*aktu&#xFFFD; (*aktu&#xFFFD; (*aktu&#xFFFD; (*aktu&#xFFFD; (*aktu&#xFFFD; (*aktu&#xFFFD; (*aktu&#xFFFD; (*aktu&#xFFFD; (*aktu&#xFFFD; (*aktu&#xFFFD; (*aktu&#xFFFD; (*aktu&#xFFFD; (*aktu&#xFFFD; (*aktu&#xFFFD; (*aktu&#xFFFD; (*aktu&#xFFFD; (*aktu&#xFFFD; (*aktu&#xFFFD; (*aktu&#xFFFD; (*aktu&#xFFFD; (*aktu&#xFFFD; (*aktu&#xFFFD; (*aktu&#xFFFD; (*aktu&#xFFFD; (*aktu&#xFFFD; (*aktu&#xFFFD; (*aktu&#xFFFD; (*aktu&#xFFFD; (*aktu&#xFFFD; (*aktu&#xFFFD; (*aktu&#xFFFD; (*aktu&#xFFFD; (*aktu&#xFFFD; (*aktu&#xFFFD; (*aktu&#xFFFD; (*aktu&#xFFFD; (*aktu&#xFFFD; (*aktu&#xFFFD; (*aktu&#xFFFD; (*aktu&#xFFFD; (*aktu&#xFFFD; (*aktu&#xFFFD; (*aktu&#xFFFD; (*aktu&#xFFFD; (*aktu&#xFFFD; (*aktu&#xFFFD; (*aktu&#xFFFD; (*aktu&#xFFFD; (*aktu&#xFFFD; (*aktu&#xFFFD; (*aktu&#xFFFD; (*aktu&#xFFFD; (*aktu&#xFFFD; (*aktu&#xFFFD; (*aktu&#xFFFD; (*aktu&#xFFFD; (*aktu&#xFFFD; (*aktu&#xFFFD; (*aktu&#xFFFD; (*aktu&#xFFFD; (*aktu&#xFFFD; (*aktu&#xFFFD; (*aktu&#xFFFD; (*aktu&#xFFFD; (*aktu&#xFFFD; (*aktu&#xFFFD; (*aktu&#xFFFD; (*aktu&#xFFFD; (*aktu&#xFFFD; (*aktu&#xFFFD; (*aktu&#xFFFD; (*aktu&#xFFFD; (*aktu&#xFFFD; (*aktu&#xFFFD; (*aktu&#xFFFD; (*aktu&#xFFFD; (*aktu&#xFFFD; (*aktu&#xFFFD; (*aktu&#xFFFD; (*aktu&#xFFFD; (*aktu&#xFFFD; (*aktu&#xFFFD; (*aktu&#xFFFD; (*aktu&#xFFFD; (*aktu&#xFFFD; (*aktu&#xFFFD; (*aktu&#xFFFD; (*aktu&#xFFFD; (*aktu&#xFFFD; (*aktu&#xFFFD; (*aktu&#xFFFD; (*aktu&#xFFFD; (*aktu&#xFFFD; (*aktu&#xFFFD; (*aktu&#xFFFD; (*aktu&#xFFFD; (*aktu&#xFFFD; (*aktu&#xFFFD; (*aktu&#xFFFD; (*aktu&#xFFFD; (*aktu&#xFFFD; (*aktu&#xFFFD; (*aktu&#xFFFD; (*aktu&#xFFFD; (*aktu&#xFFFD; (*aktu&#xFFFD; (*aktu&#xFFFD; (*aktu&#xFFFD; (*aktu&#xFFFD; (*aktu&#xFFFD; (*aktu&#xFFFD; (*aktu&#xFFFD; (*aktu&#xFFFD; (*aktu&#xFFFD; (*aktu&#xFFFD; (*aktu&#xFFFD; (*aktu&#xFFFD; (*aktu&#xFFFD; (*aktu&#xFFFD; (*aktu&#xFFFD; (*aktu&#xFFFD; (*aktu&#xFFFD; (*aktu&#xFFFD; (*aktu&#xFFFD; (*aktu&#xFFFD; (*aktu&#xFFFD; (*aktu&#xFFFD; (*aktu&#xFFFD; (*aktu&#xFFFD; (*aktu&#xFFFD; (*aktu&#xFFFD; (*aktu&#xFFFD; (*aktu&#xFFFD; (*aktu&#xFFFD; (*aktu&#xFFFD; (*aktu&#xFFFD; (*aktu&#xFFFD; (*aktu&#xFFFD; (*aktu&#xFFFD; (*aktu&#xFFFD; (*aktu&#xFFFD; (*aktu&#xFFFD; (*aktu&#xFFFD; (*aktu&#xFFFD; (*aktu&#xFFFD; (*aktu&#xFFFD; (*aktu&#xFFFD; (*aktu&#xFFFD; (*aktu&#xFFFD; (*aktu&#xFFFD; (*aktu&#xFFFD; (*aktu&#xFFFD; (*aktu&#xFFFD; (*aktu&#xFFFD; (*aktu&#xFFFD; (*aktu&#xFFFD; (*aktu&#xFFFD; (*aktu&#xFFFD; (*aktu&#xFFFD; (*aktu&#xFFFD; (*aktu&#xFFFD; (*aktu&#xFFFD; (*aktu&#xFFFD; (*aktu&#xFFFD; (*aktu&#xFFFD; (*aktu&#xFFFD; (*aktu&#xFFFD; (*aktu&#xFFFD; (*aktu&#xFFFD; (*aktu&#xFFFD; (*aktu&#xFFFD; (*aktu&#xFFFD; (*aktu&#xFFFD; (*aktu&#xFFFD; (*aktu&#xFFFD; (*aktu&#xFFFD; (*aktu&#xFFFD; (*aktu&#xFFFD; (*aktu&#xFFFD; (*aktu&#xFFFD; (*aktu&#xFFFD; (*aktu&#xFFFD; (*aktu&#xFFFD; (*aktu&#xFFFD; (*aktu&#xFFFD; (*aktu&#xFFFD; (*aktu&#xFFFD; (*aktu&#xFFFD; (*aktu&#xFFFD; (*aktu&#xFFFD; (*aktu&#xFFFD; (*aktu&#xFFFD; (*aktu&#xFFFD; (*aktu&#xFFFD; (*aktu&#xFFFD; (*aktu&#xFFFD; (*aktu&#xFFFD; (*aktu&#xFFFD; (*aktu&#xFFFD; (*aktu&#xFFFD; (*aktu&#xFFFD; (*aktu&#xFFFD; (*aktu&#xFFFD; (*aktu&#xFFFD; (*aktu&#xFFFD; (*aktu&#xFFFD; (*aktu&#xFFFD; (*aktu&#xFFFD; (*aktu&#xFFFD; (*aktu&#xFFFD; (*aktu&#xFFFD; (*aktu&#xFFFD; (*aktu&#xFFFD; (*aktu&#xFFFD; (*aktu&#xFFFD; (*aktu&#xFFFD; (*aktu&#xFFFD; (*aktu&#xFFFD; (*aktu&#xFFFD; (*aktu&#xFFFD; (*aktu&#xFFFD; (*aktu&#xFFFD; (*aktu&#xFFFD; (*aktu&#xFFFD; (*aktu&#xFFFD; (*aktu&#xFFFD; (*aktu&#xFFFD; (*aktu&#xFFFD; (*aktu&#xFFFD; (*aktu&#xFFFD; (*aktu&#xFFFD; (*aktu&#xFFFD; (*aktu&#xFFFD; (*aktu&#xFFFD; (*aktu&#xFFFD; (*aktu&#xFFFD; (*aktu&#xFFFD; (*aktu&#xFFFD; (*aktu&#xFFFD; (*aktu&#xFFFD; (*aktu&#xFFFD; (*aktu&#xFFFD; (*aktu&#xFFFD; (*aktu&#xFFFD; (*aktu&#xFFFD; (*aktu&#xFFFD; (*aktu&#xFFFD; (*aktu&#xFFFD; (*aktu&#xFFFD; (*aktu&#xFFFD; (*aktu&#xFFFD; (*aktu&#xFFFD; (*aktu&#xFFFD; (*aktu&#xFFFD; (*aktu&#xFFFD; (*aktu&#xFFFD; (*aktu&#xFFFD; (*aktu&#xFFFD; (*aktu&#xFFFD; (*aktu&#xFFFD; (*aktu&#xFFFD; (*aktu&#xFFFD; (*aktu&#xFFFD; (*aktu&#xFFFD; (*aktu&#xFFFD; (*aktu&#xFFFD; (*aktu&#xFFFD; (*aktu&#xFFFD; (*aktu&#xFFFD; (*aktu&#xFFFD; (*aktu&#xFFFD; (*aktu&#xFFFD; (*aktu&#xFFFD; (*aktu&#xFFFD; (*aktu&#xFFFD; (*aktu&#xFFFD; (*aktu&#xFFFD; (*aktu&#xFFFD; (*aktu&#xFFFD; (*aktu&#xFFFD; (*aktu&#xFFFD; (*aktu&#xFFFD; (*aktu&#xFFFD; (*aktu&#xFFFD; (*aktu&#xFFFD; (*aktu&#xFFFD; (*aktu&#xFFFD; (*aktu&#xFFFD; (*aktu&#xFFFD; (*aktu&#xFFFD; (*aktu&#xFFFD; (*aktu&#xFFFD; (*aktu&#xFFFD; (*aktu&#xFFFD; (*aktu&#xFFFD; (*aktu&#xFFFD; (*aktu&#xFFFD; (*aktu&#xFFFD; (*aktu&#xFFFD; (*aktu&#xFFFD; (*aktu&#xFFFD; (*aktu&#xFFFD; (*aktu&#xFFFD; (*aktu&#xFFFD; (*aktu&#xFFFD; (*aktu&#xFFFD; (*aktu&#xFFFD; (*aktu&#xFFFD; (*aktu&#xFFFD; (*aktu&#xFFFD; (*aktu&#xFFFD; (*aktu&#xFFFD; (*aktu&#xFFFD; (*aktu&#xFFFD; (*aktu&#xFFFD; (*aktu&#xFFFD; (*aktu&#xFFFD; (*aktu&#xFFFD; (*aktu&#xFFFD; (*aktu&#xFFFD; (*aktu&#xFFFD; (*aktu&#xFFFD; (*aktu&#xFFFD; (*aktu&#xFFFD; (*aktu&#xFFFD; (*aktu&#xFFFD; (*aktu&#xFFFD; (*aktu&#xFFFD; (*aktu&#xFFFD; (*aktu&#xFFFD; (*aktu&#xFFFD; (*aktu&#xFFFD; (*aktu&#xFFFD; (*aktu&#xFFFD; (*aktu&#xFFFD; (*aktu&#xFFFD; (*aktu&#xFFFD; (*aktu&#xFFFD; (*aktu&#xFFFD; (*aktu&#xFFFD; (*aktu&#xFFFD; (*aktu&#xFFFD; (*aktu&#xFFFD; (*aktu&#xFFFD; (*aktu&#xFFFD; (*aktu&#xFFFD; (*aktu&#xFFFD; (*aktu&#xFFFD; (*aktu&#xFFFD; (*aktu&#xFFFD; (*aktu&#xFFFD; (*aktu&#xFFFD; (*aktu&#xFFFD; (*aktu&#xFFFD; (*aktu&#xFFFD; (*aktu&#xFFFD; (*aktu&#xFFFD; (*aktu&#xFFFD; (*aktu&#xFFFD; (*aktu&#xFFFD; (*aktu&#xFFFD; (*aktu&#xFFFD; (*aktu&#xFFFD; (*aktu&#xFFFD; (*aktu&#xFFFD; (*aktu&#xFFFD; (*aktu&#xFFFD; (*aktu&#xFFFD; (*aktu&#xFFFD; (*aktu&#xFFFD; (*aktu&#xFFFD; (*aktu&#xFFFD; (*aktu&#xFFFD; (*aktu&#xFFFD; (*aktu&#xFFFD; (*aktu&#xFFFD; (*aktu&#xFFFD; (*aktu&#xFFFD; (*aktu&#xFFFD; (*aktu&#xFFFD; (*aktu&#xFFFD; (*aktu&#xFFFD; (*aktu&#xFFFD; (*aktu&#xFFFD; (*aktu&#xFFFD; (*aktu&#xFFFD; (*aktu&#xFFFD; (*aktu&#xFFFD; (*aktu&#xFFFD; (*aktu&#xFFFD; (*aktu&#xFFFD; (*aktu&#xFFFD; (*aktu&#xFFFD; (*aktu&#xFFFD; (*aktu&#xFFFD; (*aktu&#xFFFD; (*aktu&#xFFFD; (*aktu&#xFFFD; (*aktu&#xFFFD; (*aktu&#xFFFD; (*aktu&#xFFFD; (*aktu&#xFFFD; (*aktu&#xFFFD; (*aktu&#xFFFD; (*aktu&#xFFFD; (*aktu&#xFFFD; (*aktu&#xFFFD; (*aktu&#xFFFD; (*aktu&#xFFFD; (*aktu&#xFFFD; (*aktu&#xFFFD; (*aktu&#xFFFD; (*aktu&#xFFFD; (*aktu&#xFFFD; (*aktu&#xFFFD; (*aktu&#xFFFD; (*aktu&#xFFFD; (*aktu&#xFFFD; (*aktu&#xFFFD; (*aktu&#xFFFD; (*aktu&#xFFFD; (*aktu&#xFFFD; (*aktu&#xFFFD; (*aktu&#xFFFD; (*aktu&#xFFFD; (*aktu&#xFFFD; (*aktu&#xFFFD; (*aktu&#xFFFD; (*aktu&#xFFFD; (*aktu&#xFFFD; (*aktu&#xFFFD; (*aktu&#xFFFD; (*aktu&#xFFFD; (*aktu&#xFFFD; (*aktu&#xFFFD; (*aktu&#xFFFD; (*aktu&#xFFFD; (*aktu&#xFFFD; (*aktu&#xFFFD; (*aktu&#xFFFD; (*aktu&#xFFFD; (*aktu&#xFFFD; (*aktu&#xFFFD; (*aktu&#xFFFD; (*aktu&#xFFFD; (*aktu&#xFFFD; (*aktu&#xFFFD; (*aktu&#xFFFD; (*aktu&#xFFFD; (*aktu&#xFFFD; (*aktu&#xFFFD; (*aktu&#xFFFD; (*aktu&#xFFFD; (*aktu&#xFFFD; (*aktu&#xFFFD; (*aktu&#xFFFD; (*aktu&#xFFFD; (*aktu&#xFFFD; (*aktu&#xFFFD; (*aktu&#xFFFD; (*aktu&#xFFFD; (*aktu&#xFFFD; (*aktu&#xFFFD; (*aktu&#xFFFD; (*aktu&#xFFFD; (*aktu&#xFFFD; (*aktu&#xFFFD; (*aktu&#xFFFD; (*aktu&#xFFFD; (*aktu&#xFFFD; (*aktu&#xFFFD; (*aktu&#xFFFD; (*aktu&#xFFFD; (*aktu&#xFFFD; (*aktu&#xFFFD; (*aktu&#xFFFD; (*aktu&#xFFFD; (*aktu&#xFFFD; (*aktu&#xFFFD; (*aktu&#xFFFD; (*aktu&#xFFFD; (*aktu&#xFFFD; (*aktu&#xFFFD; (*aktu&#xFFFD; (*aktu&#xFFFD; (*aktu&#xFFFD; (*aktu&#xFFFD; (*aktu&#xFFFD; (*aktu&#xFFFD; (*aktu&#xFFFD; (*aktu&#xFFFD; (*aktu&#xFFFD; (*aktu&#xFFFD; (*aktu&#xFFFD; (*aktu&#xFFFD; (*aktu&#xFFFD; (*aktu&#xFFFD; (*aktu&#xFFFD; (*aktu&#xFFFD; (*aktu&#xFFFD; (*aktu&#xFFFD; (*aktu&#xFFFD; (*aktu&#xFFFD; (*aktu&#xFFFD; (*aktu&#xFFFD; (*aktu&#xFFFD; (*aktu&#xFFFD; (*aktu&#xFFFD; (*aktu&#xFFFD; (*aktu&#xFFFD; (*aktu&#xFFFD; (*aktu&#xFFFD; (*aktu&#xFFFD; (*aktu&#xFFFD; (*aktu&#xFFFD; (*aktu&#xFFFD; (*aktu&#xFFFD; (*aktu&#xFFFD; (*aktu&#xFFFD; (*aktu&#xFFFD; (*aktu&#xFFFD; (*aktu&#xFFFD; (*aktu&#xFFFD; (*aktu&#xFFFD; (*aktu&#xFFFD; (*aktu&#xFFFD; (*aktu&#xFFFD; (*aktu&#xFFFD; (*aktu&#xFFFD; (*aktu&#xFFFD; (*aktu&#xFFFD; (*aktu&#xFFFD; (*aktu&#xFFFD; (*aktu&#xFFFD; (*aktu&#xFFFD; (*aktu&#xFFFD; (*aktu&#xFFFD; (*aktu&#xFFFD; (*aktu&#xFFFD; (*aktu&#xFFFD; (*aktu&#xFFFD; (*aktu&#xFFFD; (*aktu&#xFFFD; (*aktu&#xFFFD; (*aktu&#xFFFD; (*aktu&#xFFFD; (*aktu&#xFFFD; (*aktu&#xFFFD; (*aktu&#xFFFD; (*aktu&#xFFFD; (*aktu&#xFFFD; (*aktu&#xFFFD; (*aktu&#xFFFD; (*aktu&#xFFFD; (*aktu&#xFFFD; (*aktu&#xFFFD; (*aktu&#xFFFD; (*aktu&#xFFFD; (*aktu&#xFFFD; (*aktu&#xFFFD; (*aktu&#xFFFD; (*aktu&#xFFFD; (*aktu&#xFFFD; (*aktu&#xFFFD; (*aktu&#xFFFD; (*aktu&#xFFFD; (*aktu&#xFFFD; (*aktu&#xFFFD; (*aktu&#xFFFD; (*aktu&#xFFFD; (*aktu&#xFFFD; (*aktu&#xFFFD; (*aktu&#xFFFD; (*aktu&#xFFFD; (*aktu&#xFFFD; (*aktu&#xFFFD; (*aktu&#xFFFD; (*aktu&#xFFFD; (*aktu&#xFFFD; (*aktu&#xFFFD; (*aktu&#xFFFD; (*aktu&#xFFFD; (*aktu&#xFFFD; (*aktu&#xFFFD; (*aktu&#xFFFD; (*aktu&#xFFFD; (*aktu&#xFFFD; (*aktu&#xFFFD; (*aktu&#xFFFD; (*aktu&#xFFFD; (*aktu&#xFFFD; (*aktu&#xFFFD; (*aktu&#xFFFD; (*aktu&#xFFFD; (*aktu&#xFFFD; (*aktu&#xFFFD; (*aktu&#xFFFD; (*aktu&#xFFFD; (*aktu&#xFFFD; (*aktu&#xFFFD; (*aktu&#xFFFD; (*aktu&#xFFFD; (*aktu&#xFFFD; (*aktu&#xFFFD; (*aktu&#xFFFD; (*aktu&#xFFFD; (*aktu&#xFFFD; (*aktu&#xFFFD; (*aktu&#xFFFD; (*aktu&#xFFFD; (*aktu&#xFFFD; (*aktu&#xFFFD; (*aktu&#xFFFD; (*aktu&#xFFFD; (*aktu&#xFFFD; (*aktu&#xFFFD; (*aktu&#xFFFD; (*aktu&#xFFFD; (*aktu&#xFFFD; (*aktu&#xFFFD; (*aktu&#xFFFD; (*aktu&#xFFFD; (*aktu&#xFFFD; (*aktu&#xFFFD; (*aktu&#xFFFD; (*aktu&#xFFFD; (*aktu&#xFFFD; (*aktu&#xFFFD; (*aktu&#xFFFD; (*aktu&#xFFFD; (*aktu&#xFFFD; (*aktu&#xFFFD; (*aktu&#xFFFD; (*aktu&#xFFFD; (*aktu&#xFFFD; (*aktu&#xFFFD; (*aktu&#xFFFD; (*aktu&#xFFFD; (*aktu&#xFFFD; (*aktu&#xFFFD; (*aktu&#xFFFD; (*aktu&#xFFFD; (*aktu&#xFFFD; (*aktu&#xFFFD; (*aktu&#xFFFD; (*aktu&#xFFFD; (*aktu&#xFFFD; (*aktu&#xFFFD; (*aktu&#xFFFD; (*aktu&#xFFFD; (*aktu&#xFFFD; (*aktu&#xFFFD; (*aktu&#xFFFD; (*aktu&#xFFFD; (*aktu&#xFFFD; (*aktu&#xFFFD; (*aktu&#xFFFD; (*aktu&#xFFFD; (*aktu&#xFFFD; (*aktu&#xFFFD; (*aktu&#xFFFD; (*aktu&#xFFFD; (*aktu&#xFFFD; (*aktu&#xFFFD; (*aktu&#xFFFD; (*aktu&#xFFFD; (*aktu&#xFFFD; (*aktu&#xFFFD; (*aktu&#xFFFD; (*aktu&#xFFFD; (*aktu&#xFFFD; (*aktu&#xFFFD; (*aktu&#xFFFD; (*aktu&#xFFFD; (*aktu&#xFFFD; (*aktu&#xFFFD; (*aktu&#xFFFD; (*aktu&#xFFFD; (*aktu&#xFFFD; (*aktu&#xFFFD; (*aktu&#xFFFD; (*aktu&#xFFFD; (*aktu&#xFFFD; (*aktu&#xFFFD; (*aktu&#xFFFD; (*aktu&#xFFFD; (*aktu&#xFFFD; (*aktu&#xFFFD; (*aktu&#xFFFD; (*aktu&#xFFFD; (*aktu&#xFFFD; (*aktu&#xFFFD; (*aktu&#xFFFD; (*aktu&#xFFFD; (*aktu&#xFFFD; (*aktu&#xFFFD; (*aktu&#xFFFD; (*aktu&#xFFFD; (*aktu&#xFFFD; (*aktu&#xFFFD; (*aktu&#xFFFD; (*aktu&#xFFFD; (*aktu&#xFFFD; (*aktu&#xFFFD; (*aktu&#xFFFD; (*aktu&#xFFFD; (*aktu&#xFFFD; (*aktu&#xFFFD; (*aktu&#xFFFD; (*aktu&#xFFFD; (*aktu&#xFFFD; (*aktu&#xFFFD; (*aktu&#xFFFD; (*aktu&#xFFFD; (*aktu&#xFFFD; (*aktu&#xFFFD; (*aktu&#xFFFD; (*aktu&#xFFFD; (*aktu&#xFFFD; (*aktu&#xFFFD; (*aktu&#xFFFD; (*aktu&#xFFFD; (*aktu&#xFFFD; (*aktu&#xFFFD; (*aktu&#xFFFD; (*aktu&#xFFFD; (*aktu&#xFFFD; (*aktu&#xFFFD; (*aktu&#xFFFD; (*aktu&#xFFFD; (*aktu&#xFFFD; (*aktu&#xFFFD; (*aktu&#xFFFD; (*aktu&#xFFFD; (*aktu&#xFFFD; (*aktu&#xFFFD; (*aktu&#xFFFD; (*aktu&#xFFFD; (*aktu&#xFFFD; (*aktu&#xFFFD; (*aktu&#xFFFD; (*aktu&#xFFFD; (*aktu&#xFFFD; (*aktu&#xFFFD; (*aktu&#xFFFD; (*aktu&#xFFFD; (*aktu&#xFFFD; (*aktu&#xFFFD; (*aktu&#xFFFD; (*aktu&#xFFFD; (*aktu&#xFFFD; (*aktu&#xFFFD; (*aktu&#xFFFD; (*aktu&#xFFFD; (*aktu&#xFFFD; (*aktu&#xFFFD; (*aktu&#xFFFD; (*aktu&#xFFFD; (*aktu&#xFFFD; (*aktu&#xFFFD; (*aktu&#xFFFD; (*aktu&#xFFFD; (*aktu&#xFFFD; (*aktu&#xFFFD; (*aktu&#xFFFD; (*aktu&#xFFFD; (*aktu&#xFFFD; (*aktu&#xFFFD; (*aktu&#xFFFD; (*aktu&#xFFFD; (*aktu&#xFFFD; (*aktu&#xFFFD; (*aktu&#xFFFD; (*aktu&#xFFFD; (*aktu&#xFFFD; (*aktu&#xFFFD; (*aktu&#xFFFD; (*aktu&#xFFFD; (*aktu&#xFFFD; (*aktu&#xFFFD; (*aktu&#xFFFD; (*aktu&#xFFFD; (*aktu&#xFFFD; (*aktu&#xFFFD; (*aktu&#xFFFD; (*aktu&#xFFFD; (*aktu&#xFFFD; (*aktu&#xFFFD; (*aktu&#xFFFD; (*aktu&#xFFFD; (*aktu&#xFFFD; (*aktu&#xFFFD; (*aktu&#xFFFD; (*aktu&#xFFFD; (*aktu&#xFFFD; (*aktu&#xFFFD; (*aktu&#xFFFD; (*aktu&#xFFFD; (*aktu&#xFFFD; (*aktu&#xFFFD; (*aktu&#xFFFD; (*aktu&#xFFFD; (*aktu&#xFFFD; (*aktu&#xFFFD; (*aktu&#xFFFD; (*aktu&#xFFFD; (*aktu&#xFFFD; (*aktu&#xFFFD; (*aktu&#xFFFD; (*aktu&#xFFFD; (*aktu&#xFFFD; (*aktu&#xFFFD; (*aktu&#xFFFD; (*aktu&#xFFFD; (*aktu&#xFFFD; (*aktu&#xFFFD; (*aktu&#xFFFD; (*aktu&#xFFFD; (*aktu&#xFFFD; (*aktu&#xFFFD; (*aktu&#xFFFD; (*aktu&#xFFFD; (*aktu&#xFFFD; (*aktu&#xFFFD; (*aktu&#xFFFD; (*aktu&#xFFFD; (*aktu&#xFFFD; (*aktu&#xFFFD; (*aktu&#xFFFD; (*aktu&#xFFFD; (*aktu&#xFFFD; (*aktu&#xFFFD; (*aktu&#xFFFD; (*aktu&#xFFFD; (*aktu&#xFFFD; (*aktu&#xFFFD; (*aktu&#xFFFD; (*aktu&#xFFFD; (*aktu&#xFFFD; (*aktu&#xFFFD; (*aktu&#xFFFD; (*aktu&#xFFFD; (*aktu&#xFFFD; (*aktu&#xFFFD; (*aktu&#xFFFD; (*aktu&#xFFFD; (*aktu&#xFFFD; (*aktu&#xFFFD; (*aktu&#xFFFD; (*aktu&#xFFFD; (*aktu&#xFFFD; (*aktu&#xFFFD; (*aktu&#xFFFD; (*aktu&#xFFFD; (*aktu&#xFFFD; (*aktu&#xFFFD; (*aktu&#xFFFD; (*aktu&#xFFFD; (*aktu&#xFFFD; (*aktu&#xFFFD; (*aktu&#xFFFD; (*aktu&#xFFFD; (*aktu&#xFFFD; (*aktu&#xFFFD; (*aktu&#xFFFD; (*aktu&#xFFFD; (*aktu&#xFFFD; (*aktu&#xFFFD; (*aktu&#xFFFD; (*aktu&#xFFFD; (*aktu&#xFFFD; (*aktu&#xFFFD; (*aktu&#xFFFD; (*aktu&#xFFFD; (*aktu&#xFFFD; (*aktu&#xFFFD; (*aktu&#xFFFD; (*aktu&#xFFFD; (*aktu&#xFFFD; (*aktu&#xFFFD; (*aktu&#xFFFD; (*aktu&#xFFFD; (*aktu&#xFFFD; (*aktu&#xFFFD; (*aktu&#xFFFD; (*aktu&#xFFFD; (*aktu&#xFFFD; (*aktu&#xFFFD; (*aktu&#xFFFD; (*aktu&#xFFFD; (*aktu&#xFFFD; (*aktu&#xFFFD; (*aktu&#xFFFD; (*aktu&#xFFFD; (*aktu&#xFFFD; (*aktu&#xFFFD; (*aktu&#xFFFD; (*aktu&#xFFFD; (*aktu&#xFFFD; (*aktu&#xFFFD; (*aktu&#xFFFD; (*aktu&#xFFFD; (*aktu&#xFFFD; (*aktu&#xFFFD; (*aktu&#xFFFD; (*aktu&#xFFFD; (*aktu&#xFFFD; (*aktu&#xFFFD; (*aktu&#xFFFD; (*aktu&#xFFFD; (*aktu&#xFFFD; (*aktu&#xFFFD; (*aktu&#xFFFD; (*aktu&#xFFFD; (*aktu&#xFFFD; (*aktu&#xFFFD; (*aktu&#xFFFD; (*aktu&#xFFFD; (*aktu&#xFFFD; (*aktu&#xFFFD; (*aktu&#xFFFD; (*aktu&#xFFFD; (*aktu&#xFFFD; (*aktu&#xFFFD; (*aktu&#xFFFD; (*aktu&#xFFFD; (*aktu&#xFFFD; (*aktu&#xFFFD; (*aktu&#xFFFD; (*aktu&#xFFFD; (*aktu&#xFFFD; (*aktu&#xFFFD; (*aktu&#xFFFD; (*aktu&#xFFFD; (*aktu&#xFFFD; (*aktu&#xFFFD; (*aktu&#xFFFD; (*aktu&#xFFFD; (*aktu&#xFFFD; (*aktu&#xFFFD; (*aktu&#xFFFD; (*aktu&#xFFFD; (*aktu&#xFFFD; (*aktu&#xFFFD; (*aktu&#xFFFD; (*aktu&#xFFFD; (*aktu&#xFFFD; (*aktu&#xFFFD; (*aktu&#xFFFD; (*aktu&#xFFFD; (*aktu&#xFFFD; (*aktu&#xFFFD; (*aktu&#xFFFD; (*aktu&#xFFFD; (*aktu&#xFFFD; (*aktu&#xFFFD; (*aktu&#xFFFD; (*aktu&#xFFFD; (*aktu&#xFFFD; (*aktu&#xFFFD; (*aktu&#xFFFD; (*aktu&#xFFFD; (*aktu&#xFFFD; (*aktu&#xFFFD; (*aktu&#xFFFD; (*aktu&#xFFFD; (*aktu&#xFFFD; (*aktu&#xFFFD; (*aktu&#xFFFD; (*aktu&#xFFFD; (*aktu&#xFFFD; (*aktu&#xFFFD; (*aktu&#xFFFD; (*aktu&#xFFFD; (*aktu&#xFFFD; (*aktu&#xFFFD; (*aktu&#xFFFD; (*aktu&#xFFFD; (*aktu&#xFFFD; (*aktu&#xFFFD; (*aktu&#xFFFD; (*aktu&#xFFFD; (*aktu&#xFFFD; (*aktu&#xFFFD; (*aktu&#xFFFD; (*aktu&#xFFFD; (*aktu&#xFFFD; (*aktu&#xFFFD; (*aktu&#xFFFD; (*aktu&#xFFFD; (*aktu&#xFFFD; (*aktu&#xFFFD; (*aktu&#xFFFD; (*aktu&#xFFFD; (*aktu&#xFFFD; (*aktu&#xFFFD; (*aktu&#xFFFD; (*aktu&#xFFFD; (*aktu&#xFFFD; (*aktu&#xFFFD; (*aktu&#xFFFD; (*aktu&#xFFFD; (*aktu&#xFFFD; (*aktu&#xFFFD; (*aktu&#xFFFD; (*aktu&#xFFFD; (*aktu&#xFFFD; (*aktu&#xFFFD; (*aktu&#xFFFD; (*aktu&#xFFFD; (*aktu&#xFFFD; (*aktu&#xFFFD; (*aktu&#xFFFD; (*aktu&#xFFFD; (*aktu&#xFFFD; (*aktu&#xFFFD; (*aktu&#xFFFD; (*aktu&#xFFFD; (*aktu&#xFFFD; (*aktu&#xFFFD; (*aktu&#xFFFD; (*aktu&#xFFFD; (*aktu&#xFFFD; (*aktu&#xFFFD; (*aktu&#xFFFD; (*aktu&#xFFFD; (*aktu&#xFFFD; (*aktu&#xFFFD; (*aktu&#xFFFD; (*aktu&#xFFFD; (*aktu&#xFFFD; (*aktu&#xFFFD; (*aktu&#xFFFD; (*aktu&#xFFFD; (*aktu&#xFFFD; (*aktu&#xFFFD; (*aktu&#xFFFD; (*aktu&#xFFFD; (*aktu&#xFFFD; (*aktu&#xFFFD; (*aktu&#xFFFD; (*aktu&#xFFFD; (*aktu&#xFFFD; (*aktu&#xFFFD; (*aktu&#xFFFD; (*aktu&#xFFFD; (*aktu&#xFFFD; (*aktu&#xFFFD; (*aktu&#xFFFD; (*aktu&#xFFFD; (*aktu&#xFFFD; (*aktu&#xFFFD; (*aktu&#xFFFD; (*aktu&#xFFFD; (*aktu&#xFFFD; (*aktu&#xFFFD; (*aktu&#xFFFD; (*aktu&#xFFFD; (*aktu&#xFFFD; (*aktu&#xFFFD; (*aktu&#xFFFD; (*aktu&#xFFFD; (*aktu&#xFFFD; (*aktu&#xFFFD; (*aktu&#xFFFD; (*aktu&#xFFFD; (*aktu&#xFFFD; (*aktu&#xFFFD; (*aktu&#xFFFD; (*aktu&#xFFFD; (*aktu&#xFFFD; (*aktu&#xFFFD; (*aktu&#xFFFD; (*aktu&#xFFFD; (*aktu&#xFFFD; (*aktu&#xFFFD; (*aktu&#xFFFD; (*aktu&#xFFFD; (*aktu&#xFFFD; (*aktu&#xFFFD; (*aktu&#xFFFD; (*aktu&#xFFFD; (*aktu&#xFFFD; (*aktu&#xFFFD; (*aktu&#xFFFD; (*aktu&#xFFFD; (*aktu&#xFFFD; (*aktu&#xFFFD; (*aktu&#xFFFD; (*aktu&#xFFFD; (*aktu&#xFFFD; (*aktu&#xFFFD; (*aktu&#xFFFD; (*aktu&#xFFFD; (*aktu&#xFFFD; (*aktu&#xFFFD; (*aktu&#xFFFD; (*aktu&#xFFFD; (*aktu&#xFFFD; (*aktu&#xFFFD; (*aktu&#xFFFD; (*aktu&#xFFFD; (*aktu&#xFFFD; (*aktu&#xFFFD; (*aktu&#xFFFD; (*aktu&#xFFFD; (*aktu&#xFFFD; (*aktu&#xFFFD; (*aktu&#xFFFD; (*aktu&#xFFFD; (*aktu&#xFFFD; (*aktu&#xFFFD; (*aktu&#xFFFD; (*aktu&#xFFFD; (*aktu&#xFFFD; (*aktu&#xFFFD; (*aktu&#xFFFD; (*aktu&#xFFFD; (*aktu&#xFFFD; (*aktu&#xFFFD; (*aktu&#xFFFD; (*aktu&#xFFFD; (*aktu&#xFFFD; (*aktu&#xFFFD; (*aktu&#xFFFD; (*aktu&#xFFFD; (*aktu&#xFFFD; (*aktu&#xFFFD; (*aktu&#xFFFD; (*aktu&#xFFFD; (*aktu&#xFFFD; (*aktu&#xFFFD; (*aktu&#xFFFD; (*aktu&#xFFFD; (*aktu&#xFFFD; (*aktu&#xFFFD; (*aktu&#xFFFD; (*aktu&#xFFFD; (*aktu&#xFFFD; (*aktu&#xFFFD; (*aktu&#xFFFD; (*aktu&#xFFFD; (*aktu&#xFFFD; (*aktu&#xFFFD; (*aktu&#xFFFD; (*aktu&#xFFFD; (*aktu&#xFFFD; (*aktu&#xFFFD; (*aktu&#xFFFD; (*aktu&#xFFFD; (*aktu&#xFFFD; (*aktu&#xFFFD; (*aktu&#xFFFD; (*aktu&#xFFFD; (*aktu&#xFFFD; (*aktu&#xFFFD; (*aktu&#xFFFD; (*aktu&#xFFFD; (*aktu&#xFFFD; (*aktu&#xFFFD; (*aktu&#xFFFD; (*aktu&#xFFFD; (*aktu&#xFFFD; (*aktu&#xFFFD; (*aktu&#xFFFD; (*aktu&#xFFFD; (*aktu&#xFFFD; (*aktu&#xFFFD; (*aktu&#xFFFD; (*aktu&#xFFFD; (*aktu&#xFFFD; (*aktu&#xFFFD; (*aktu&#xFFFD; (*aktu&#xFFFD; (*aktu&#xFFFD; (*aktu&#xFFFD; (*aktu&#xFFFD; (*aktu&#xFFFD; (*aktu&#xFFFD; (*aktu&#xFFFD; (*aktu&#xFFFD; (*aktu&#xFFFD; (*aktu&#xFFFD; (*aktu&#xFFFD; (*aktu&#xFFFD; (*aktu&#xFFFD; (*aktu&#xFFFD; (*aktu&#xFFFD; (*aktu&#xFFFD; (*aktu&#xFFFD; (*aktu&#xFFFD; (*aktu&#xFFFD; (*aktu&#xFFFD; (*aktu&#xFFFD; (*aktu&#xFFFD; (*aktu&#xFFFD; (*aktu&#xFFFD; (*aktu&#xFFFD; (*aktu&#xFFFD; (*aktu&#xFFFD; (*aktu&#xFFFD; (*aktu&#xFFFD; (*aktu&#xFFFD; (*aktu&#xFFFD; (*aktu&#xFFFD; (*aktu&#xFFFD; (*aktu&#xFFFD; (*aktu&#xFFFD; (*aktu&#xFFFD; (*aktu&#xFFFD; (*aktu&#xFFFD; (*aktu&#xFFFD; (*aktu&#xFFFD; (*aktu&#xFFFD; (*aktu&#xFFFD; (*aktu&#xFFFD; (*aktu&#xFFFD; (*aktu&#xFFFD; (*aktu&#xFFFD; (*aktu&#xFFFD; (*aktu&#xFFFD; (*aktu&#xFFFD; (*aktu&#xFFFD; (*aktu&#xFFFD; (*aktu&#xFFFD; (*aktu&#xFFFD; (*aktu&#xFFFD; (*aktu&#xFFFD; (*aktu&#xFFFD; (*aktu&#xFFFD; (*aktu&#xFFFD; (*aktu&#xFFFD; (*aktu&#xFFFD; (*aktu&#xFFFD; (*aktu&#xFFFD; (*aktu&#xFFFD; (*aktu&#xFFFD; (*aktu&#xFFFD; (*aktu&#xFFFD; (*aktu&#xFFFD; (*aktu&#xFFFD; (*aktu&#xFFFD; (*aktu&#xFFFD; (*aktu&#xFFFD; (*aktu&#xFFFD; (*aktu&#xFFFD; (*aktu&#xFFFD; (*aktu&#xFFFD; (*aktu&#xFFFD; (*aktu&#xFFFD; (*aktu&#xFFFD; (*aktu&#xFFFD; (*aktu&#xFFFD; (*aktu&#xFFFD; (*aktu&#xFFFD; (*aktu&#xFFFD; (*aktu&#xFFFD; (*aktu&#xFFFD; (*aktu&#xFFFD; (*aktu&#xFFFD; (*aktu&#xFFFD; (*aktu&#xFFFD; (*aktu&#xFFFD; (*aktu&#xFFFD; (*aktu&#xFFFD; (*aktu&#xFFFD; (*aktu&#xFFFD; (*aktu&#xFFFD; (*aktu&#xFFFD; (*aktu&#xFFFD; (*aktu&#xFFFD; (*aktu&#xFFFD; (*aktu&#xFFFD; (*aktu&#xFFFD; (*aktu&#xFFFD; (*aktu&#xFFFD; (*aktu&#xFFFD; (*aktu&#xFFFD; (*aktu&#xFFFD; (*aktu&#xFFFD; (*aktu&#xFFFD; (*aktu&#xFFFD; (*aktu&#xFFFD; (*aktu&#xFFFD; (*aktu&#xFFFD; (*aktu&#xFFFD; (*aktu&#xFFFD; (*aktu&#xFFFD; (*aktu&#xFFFD; (*aktu&#xFFFD; (*aktu&#xFFFD; (*aktu&#xFFFD; (*aktu&#xFFFD; (*aktu&#xFFFD; (*aktu&#xFFFD; (*aktu&#xFFFD; (*aktu&#xFFFD; (*aktu&#xFFFD; (*aktu&#xFFFD; (*aktu&#xFFFD; (*aktu&#xFFFD; (*aktu&#xFFFD; (*aktu&#xFFFD; (*aktu&#xFFFD; (*aktu&#xFFFD; (*aktu&#xFFFD; (*aktu&#xFFFD; (*aktu&#xFFFD; (*aktu&#xFFFD; (*aktu&#xFFFD; (*aktu&#xFFFD; (*aktu&#xFFFD; (*aktu&#xFFFD; (*aktu&#xFFFD; (*aktu&#xFFFD; (*aktu&#xFFFD; (*aktu&#xFFFD; (*aktu&#xFFFD; (*aktu&#xFFFD; (*aktu&#xFFFD; (*aktu&#xFFFD; (*aktu&#xFFFD; (*aktu&#xFFFD; (*aktu&#xFFFD; (*aktu&#xFFFD; (*aktu&#xFFFD; (*aktu&#xFFFD; (*aktu&#xFFFD; (*aktu&#xFFFD; (*aktu&#xFFFD; (*aktu&#xFFFD; (*aktu&#xFFFD; (*aktu&#xFFFD; (*aktu&#xFFFD; (*aktu&#xFFFD; (*aktu&#xFFFD; (*aktu&#xFFFD; (*aktu&#xFFFD; (*aktu&#xFFFD; (*aktu&#xFFFD; (*aktu&#xFFFD; (*aktu&#xFFFD; (*aktu&#xFFFD; (*aktu&#xFFFD; (*aktu&#xFFFD; (*aktu&#xFFFD; (*aktu&#xFFFD; (*aktu&#xFFFD; (*aktu&#xFFFD; (*aktu&#xFFFD; (*aktu&#xFFFD; (*aktu&#xFFFD; (*aktu&#xFFFD; (*aktu&#xFFFD; (*aktu&#xFFFD; (*aktu&#xFFFD; (*aktu&#xFFFD; (*aktu&#xFFFD; (*aktu&#xFFFD; (*aktu&#xFFFD; (*aktu&#xFFFD; (*aktu&#xFFFD; (*aktu&#xFFFD; (*aktu&#xFFFD; (*aktu&#xFFFD; (*aktu&#xFFFD; (*aktu&#xFFFD; (*aktu&#xFFFD; (*aktu&#xFFFD; (*aktu&#xFFFD; (*aktu&#xFFFD; (*aktu&#xFFFD; (*aktu&#xFFFD; (*aktu&#xFFFD; (*aktu&#xFFFD; (*aktu&#xFFFD; (*aktu&#xFFFD; (*aktu&#xFFFD; (*aktu&#xFFFD; (*aktu&#xFFFD; (*aktu&#xFFFD; (*aktu&#xFFFD; (*aktu&#xFFFD; (*aktu&#xFFFD; (*aktu&#xFFFD; (*aktu&#xFFFD; (*aktu&#xFFFD; (*aktu&#xFFFD; (*aktu&#xFFFD; (*aktu&#xFFFD; (*aktu&#xFFFD; (*aktu&#xFFFD; (*aktu&#xFFFD; (*aktu&#xFFFD; (*aktu&#xFFFD; (*aktu&#xFFFD; (*aktu&#xFFFD; (*aktu&#xFFFD; (*aktu&#xFFFD; (*aktu&#xFFFD; (*aktu&#xFFFD; (*aktu&#xFFFD; (*aktu&#xFFFD; (*aktu&#xFFFD; (*aktu&#xFFFD; (*aktu&#xFFFD; (*aktu&#xFFFD; (*aktu&#xFFFD; (*aktu&#xFFFD; (*aktu&#xFFFD; (*aktu&#xFFFD; (*aktu&#xFFFD; (*aktu&#xFFFD; (*aktu&#xFFFD; (*aktu&#xFFFD; (*aktu&#xFFFD; (*aktu&#xFFFD; (*aktu&#xFFFD; (*aktu&#xFFFD; (*aktu&#xFFFD; (*aktu&#xFFFD; (*aktu&#xFFFD; (*aktu&#xFFFD; (*aktu&#xFFFD; (*aktu&#xFFFD; (*aktu&#xFFFD; (*aktu&#xFFFD; (*aktu&#xFFFD; (*aktu&#xFFFD; (*aktu&#xFFFD; (*aktu&#xFFFD; (*aktu&#xFFFD; (*aktu&#xFFFD; (*aktu&#xFFFD; (*aktu&#xFFFD; (*aktu&#xFFFD; (*aktu&#xFFFD; (*aktu&#xFFFD; (*aktu&#xFFFD; (*aktu&#xFFFD; (*aktu&#xFFFD; (*aktu&#xFFFD; (*aktu&#xFFFD; (*aktu&#xFFFD; (*aktu&#xFFFD; (*aktu&#xFFFD; (*aktu&#xFFFD; (*aktu&#xFFFD; (*aktu&#xFFFD; (*aktu&#xFFFD; (*aktu&#xFFFD; (*aktu&#xFFFD; (*aktu&#xFFFD; (*aktu&#xFFFD; (*aktu&#xFFFD; (*aktu&#xFFFD; (*aktu&#xFFFD; (*aktu&#xFFFD; (*aktu&#xFFFD; (*aktu&#xFFFD; (*aktu&#xFFFD; (*aktu&#xFFFD; (*aktu&#xFFFD; (*aktu&#xFFFD; (*aktu&#xFFFD; (*aktu&#xFFFD; (*aktu&#xFFFD; (*aktu&#xFFFD; (*aktu&#xFFFD; (*aktu&#xFFFD; (*aktu&#xFFFD; (*aktu&#xFFFD; (*aktu&#xFFFD; (*aktu&#xFFFD; (*aktu&#xFFFD; (*aktu&#xFFFD; (*aktu&#xFFFD; (*aktu&#xFFFD; (*aktu&#xFFFD; (*aktu&#xFFFD; (*aktu&#xFFFD; (*aktu&#xFFFD; (*aktu&#xFFFD; (*aktu&#xFFFD; (*aktu&#xFFFD; (*aktu&#xFFFD; (*aktu&#xFFFD; (*aktu&#xFFFD; (*aktu&#xFFFD; (*aktu&#xFFFD; (*aktu&#xFFFD; (*aktu&#xFFFD; (*aktu&#xFFFD; (*aktu&#xFFFD; (*aktu&#xFFFD; (*aktu&#xFFFD; (*aktu&#xFFFD; (*aktu&#xFFFD; (*aktu&#xFFFD; (*aktu&#xFFFD; (*aktu&#xFFFD; (*aktu&#xFFFD; (*aktu&#xFFFD; (*aktu&#xFFFD; (*aktu&#xFFFD; (*aktu&#xFFFD; (*aktu&#xFFFD; (*aktu&#xFFFD; (*aktu&#xFFFD; (*aktu&#xFFFD; (*aktu&#xFFFD; (*aktu&#xFFFD; (*aktu&#xFFFD; (*aktu&#xFFFD; (*aktu&#xFFFD; (*aktu&#xFFFD; (*aktu&#xFFFD; (*aktu&#xFFFD; (*aktu&#xFFFD; (*aktu&#xFFFD; (*aktu&#xFFFD; (*aktu&#xFFFD; (*aktu&#xFFFD; (*aktu&#xFFFD; (*aktu&#xFFFD; (*aktu&#xFFFD; (*aktu&#xFFFD; (*aktu&#xFFFD; (*aktu&#xFFFD; (*aktu&#xFFFD; (*aktu&#xFFFD; (*aktu&#xFFFD; (*aktu&#xFFFD; (*aktu&#xFFFD; (*aktu&#xFFFD; (*aktu&#xFFFD; (*aktu&#xFFFD; (*aktu&#xFFFD; (*aktu&#xFFFD; (*aktu&#xFFFD; (*aktu&#xFFFD; (*aktu&#xFFFD; (*aktu&#xFFFD; (*aktu&#xFFFD; (*aktu&#xFFFD; (*aktu&#xFFFD; (*aktu&#xFFFD; (*aktu&#xFFFD; (*aktu&#xFFFD; (*aktu&#xFFFD; (*aktu&#xFFFD; (*aktu&#xFFFD; (*aktu&#xFFFD; (*aktu&#xFFFD; (*aktu&#xFFFD; (*aktu&#xFFFD; (*aktu&#xFFFD; (*aktu&#xFFFD; (*aktu&#xFFFD; (*aktu&#xFFFD; (*aktu&#xFFFD; (*aktu&#xFFFD; (*aktu&#xFFFD; (*aktu&#xFFFD; (*aktu&#xFFFD; (*aktu&#xFFFD; (*aktu&#xFFFD; (*aktu&#xFFFD; (*aktu&#xFFFD; (*aktu&#xFFFD; (*aktu&#xFFFD; (*aktu&#xFFFD; (*aktu&#xFFFD; (*aktu&#xFFFD; (*aktu&#xFFFD; (*aktu&#xFFFD; (*aktu&#xFFFD; (*aktu&#xFFFD; (*aktu&#xFFFD; (*aktu&#xFFFD; (*aktu&#xFFFD; (*aktu&#xFFFD; (*aktu&#xFFFD; (*aktu&#xFFFD; (*aktu&#xFFFD; (*aktu&#xFFFD; (*aktu&#xFFFD; (*aktu&#xFFFD; (*aktu&#xFFFD; (*aktu&#xFFFD; (*aktu&#xFFFD; (*aktu&#xFFFD; (*aktu&#xFFFD; (*aktu&#xFFFD; (*aktu&#xFFFD; (*aktu&#xFFFD; (*aktu&#xFFFD; (*aktu&#xFFFD; (*aktu&#xFFFD; (*aktu&#xFFFD; (*aktu&#xFFFD; (*aktu&#xFFFD; (*aktu&#xFFFD; (*aktu&#xFFFD; (*aktu&#xFFFD; (*aktu&#xFFFD; (*aktu&#xFFFD; (*aktu&#xFFFD; (*aktu&#xFFFD; (*aktu&#xFFFD; (*aktu&#xFFFD; (*aktu&#xFFFD; (*aktu&#xFFFD; (*aktu&#xFFFD; (*aktu&#xFFFD; (*aktu&#xFFFD; (*aktu&#xFFFD; (*aktu&#xFFFD; (*aktu&#xFFFD; (*aktu&#xFFFD; (*aktu&#xFFFD; (*aktu&#xFFFD; (*aktu&#xFFFD; (*aktu&#xFFFD; (*aktu&#xFFFD; (*aktu&#xFFFD; (*aktu&#xFFFD; (*aktu&#xFFFD; (*aktu&#xFFFD; (*aktu&#xFFFD; (*aktu&#xFFFD; (*aktu&#xFFFD; (*aktu&#xFFFD; (*aktu&#xFFFD; (*aktu&#xFFFD; (*aktu&#xFFFD; (*aktu&#xFFFD; (*aktu&#xFFFD; (*aktu&#xFFFD; (*aktu&#xFFFD; (*aktu&#xFFFD; (*aktu&#xFFFD; (*aktu&#xFFFD; (*aktu&#xFFFD; (*aktu&#xFFFD; (*aktu&#xFFFD; (*aktu&#xFFFD; (*aktu&#xFFFD; (*aktu&#xFFFD; (*aktu&#xFFFD; (*aktu&#xFFFD; (*aktu&#xFFFD; (*aktu&#xFFFD; (*aktu&#xFFFD; (*aktu&#xFFFD; (*aktu&#xFFFD; (*aktu&#xFFFD; (*aktu&#xFFFD; (*aktu&#xFFFD; (*aktu&#xFFFD; (*aktu&#xFFFD; (*aktu&#xFFFD; (*aktu&#xFFFD; (*aktu&#xFFFD; (*aktu&#xFFFD; (*aktu&#xFFFD; (*aktu&#xFFFD; (*aktu&#xFFFD; (*aktu&#xFFFD; (*aktu&#xFFFD; (*aktu&#xFFFD; (*aktu&#xFFFD; (*aktu&#xFFFD; (*aktu&#xFFFD; (*aktu&#xFFFD; (*aktu&#xFFFD; (*aktu&#xFFFD; (*aktu&#xFFFD; (*aktu&#xFFFD; (*aktu&#xFFFD; (*aktu&#xFFFD; (*aktu&#xFFFD; (*aktu&#xFFFD; (*aktu&#xFFFD; (*aktu&#xFFFD; (*aktu&#xFFFD; (*aktu&#xFFFD; (*aktu&#xFFFD; (*aktu&#xFFFD; (*aktu&#xFFFD; (*aktu&#xFFFD; (*aktu&#xFFFD; (*aktu&#xFFFD; (*aktu&#xFFFD; (*aktu&#xFFFD; (*aktu&#xFFFD; (*aktu&#xFFFD; (*aktu&#xFFFD; (*aktu&#xFFFD; (*aktu&#xFFFD; (*aktu&#xFFFD; (*aktu&#xFFFD; (*aktu&#xFFFD; (*aktu&#xFFFD; (*aktu&#xFFFD; (*aktu&#xFFFD; (*aktu&#xFFFD; (*aktu&#xFFFD; (*aktu&#xFFFD; (*aktu&#xFFFD; (*aktu&#xFFFD; (*aktu&#xFFFD; (*aktu&#xFFFD; (*aktu&#xFFFD; (*aktu&#xFFFD; (*aktu&#xFFFD; (*aktu&#xFFFD; (*aktu&#xFFFD; (*aktu&#xFFFD; (*aktu&#xFFFD; (*aktu&#xFFFD; (*aktu&#xFFFD; (*aktu&#xFFFD; (*aktu&#xFFFD; (*aktu&#xFFFD; (*aktu&#xFFFD; (*aktu&#xFFFD; (*aktu&#xFFFD; (*aktu&#xFFFD; (*aktu&#xFFFD; (*aktu&#xFFFD; (*aktu&#xFFFD; (*aktu&#xFFFD; (*aktu&#xFFFD; (*aktu&#xFFFD; (*aktu&#xFFFD; (*aktu&#xFFFD; (*aktu&#xFFFD; (*aktu&#xFFFD; (*aktu&#xFFFD; (*aktu&#xFFFD; (*aktu&#xFFFD; (*aktu&#xFFFD; (*aktu&#xFFFD; (*aktu&#xFFFD; (*aktu&#xFFFD; (*aktu&#xFFFD; (*aktu&#xFFFD; (*aktu&#xFFFD; (*aktu&#xFFFD; (*aktu&#xFFFD; (*aktu&#xFFFD; (*aktu&#xFFFD; (*aktu&#xFFFD; (*aktu&#xFFFD; (*aktu&#xFFFD; (*aktu&#xFFFD; (*aktu&#xFFFD; (*aktu&#xFFFD; (*aktu&#xFFFD; (*aktu&#xFFFD; (*aktu&#xFFFD; (*aktu&#xFFFD; (*aktu&#xFFFD; (*aktu&#xFFFD; (*aktu&#xFFFD; (*aktu&#xFFFD; (*aktu&#xFFFD; (*aktu&#xFFFD; (*aktu&#xFFFD; (*aktu&#xFFFD; (*aktu&#xFFFD; (*aktu&#xFFFD; (*aktu&#xFFFD; (*aktu&#xFFFD; (*aktu&#xFFFD; (*aktu&#xFFFD; (*aktu&#xFFFD; (*aktu&#xFFFD; (*aktu&#xFFFD; (*aktu&#xFFFD; (*aktu&#xFFFD; (*aktu&#xFFFD; (*aktu&#xFFFD; (*aktu&#xFFFD; (*aktu&#xFFFD; (*aktu&#xFFFD; (*aktu&#xFFFD; (*aktu&#xFFFD; (*aktu&#xFFFD; (*aktu&#xFFFD; (*aktu&#xFFFD; (*aktu&#xFFFD; (*aktu&#xFFFD; (*aktu&#xFFFD; (*aktu&#xFFFD; (*aktu&#xFFFD; (*aktu&#xFFFD; (*aktu&#xFFFD; (*aktu&#xFFFD; (*aktu&#xFFFD; (*aktu&#xFFFD; (*aktu&#xFFFD; (*aktu&#xFFFD; (*aktu&#xFFFD; (*aktu&#xFFFD; (*aktu&#xFFFD; (*aktu&#xFFFD; (*aktu&#xFFFD; (*aktu&#xFFFD; (*aktu&#xFFFD; (*aktu&#xFFFD; (*aktu&#xFFFD; (*aktu&#xFFFD; (*aktu&#xFFFD; (*aktu&#xFFFD; (*aktu&#xFFFD; (*aktu&#xFFFD; (*aktu&#xFFFD; (*aktu&#xFFFD; (*aktu&#xFFFD; (*aktu&#xFFFD; (*aktu&#xFFFD; (*aktu&#xFFFD; (*aktu&#xFFFD; (*aktu&#xFFFD; (*aktu&#xFFFD; (*aktu&#xFFFD; (*aktu&#xFFFD; (*aktu&#xFFFD; (*aktu&#xFFFD; (*aktu&#xFFFD; (*aktu&#xFFFD; (*aktu&#xFFFD; (*aktu&#xFFFD; (*aktu&#xFFFD; (*aktu&#xFFFD; (*aktu&#xFFFD; (*aktu&#xFFFD; (*aktu&#xFFFD; (*aktu&#xFFFD; (*aktu&#xFFFD; (*aktu&#xFFFD; (*aktu&#xFFFD; (*aktu&#xFFFD; (*aktu&#xFFFD; (*aktu&#xFFFD; (*aktu&#xFFFD; (*aktu&#xFFFD; (*aktu&#xFFFD; (*aktu&#xFFFD; (*aktu&#xFFFD; (*aktu&#xFFFD; (*aktu&#xFFFD; (*aktu&#xFFFD; (*aktu&#xFFFD; (*aktu&#xFFFD; (*aktu&#xFFFD; (*aktu&#xFFFD; (*aktu&#xFFFD; (*aktu&#xFFFD; (*aktu&#xFFFD; (*aktu&#xFFFD; (*aktu&#xFFFD; (*aktu&#xFFFD; (*aktu&#xFFFD; (*aktu&#xFFFD; (*aktu&#xFFFD; (*aktu&#xFFFD; (*aktu&#xFFFD; (*aktu&#xFFFD; (*aktu&#xFFFD; (*aktu&#xFFFD; (*aktu&#xFFFD; (*aktu&#xFFFD; (*aktu&#xFFFD; (*aktu&#xFFFD; (*aktu&#xFFFD; (*aktu&#xFFFD; (*aktu&#xFFFD; (*aktu&#xFFFD; (*aktu&#xFFFD; (*aktu&#xFFFD; (*aktu&#xFFFD; (*aktu&#xFFFD; (*aktu&#xFFFD; (*aktu&#xFFFD; (*aktu&#xFFFD; (*aktu&#xFFFD; (*aktu&#xFFFD; (*aktu&#xFFFD; (*aktu&#xFFFD; (*aktu&#xFFFD; (*aktu&#xFFFD; (*aktu&#xFFFD; (*aktu&#xFFFD; (*aktu&#xFFFD; (*aktu&#xFFFD; (*aktu&#xFFFD; (*aktu&#xFFFD; (*aktu&#xFFFD; (*aktu&#xFFFD; (*aktu&#xFFFD; (*aktu&#xFFFD; (*aktu&#xFFFD; (*aktu&#xFFFD; (*aktu&#xFFFD; (*aktu&#xFFFD; (*aktu&#xFFFD; (*aktu&#xFFFD; (*aktu&#xFFFD; (*aktu&#xFFFD; (*aktu&#xFFFD; (*aktu&#xFFFD; (*aktu&#xFFFD; (*aktu&#xFFFD; (*aktu&#xFFFD; (*aktu&#xFFFD; (*aktu&#xFFFD; (*aktu&#xFFFD; (*aktu&#xFFFD; (*aktu&#xFFFD; (*aktu&#xFFFD; (*aktu&#xFFFD; (*aktu&#xFFFD; (*aktu&#xFFFD; (*aktu&#xFFFD; (*aktu&#xFFFD; (*aktu&#xFFFD; (*aktu&#xFFFD; (*aktu&#xFFFD; (*aktu&#xFFFD; (*aktu&#xFFFD; (*aktu&#xFFFD; (*aktu&#xFFFD; (*aktu&#xFFFD; (*aktu&#xFFFD; (*aktu&#xFFFD; (*aktu&#xFFFD; (*aktu&#xFFFD; (*aktu&#xFFFD; (*aktu&#xFFFD; (*aktu&#xFFFD; (*aktu&#xFFFD; (*aktu&#xFFFD; (*aktu&#xFFFD; (*aktu&#xFFFD; (*aktu&#xFFFD; (*aktu&#xFFFD; (*aktu&#xFFFD; (*aktu&#xFFFD; (*aktu&#xFFFD; (*aktu&#xFFFD; (*aktu&#xFFFD; (*aktu&#xFFFD; (*aktu&#xFFFD; (*aktu&#xFFFD; (*aktu&#xFFFD; (*aktu&#xFFFD; (*aktu&#xFFFD; (*aktu&#xFFFD; (*aktu&#xFFFD; (*aktu&#xFFFD; (*aktu&#xFFFD; (*aktu&#xFFFD; (*aktu&#xFFFD; (*aktu&#xFFFD; (*aktu&#xFFFD; (*aktu&#xFFFD; (*aktu&#xFFFD; (*aktu&#xFFFD; (*aktu&#xFFFD; (*aktu&#xFFFD; (*aktu&#xFFFD; (*aktu&#xFFFD; (*aktu&#xFFFD; (*aktu&#xFFFD; (*aktu&#xFFFD; (*aktu&#xFFFD; (*aktu&#xFFFD; (*aktu&#xFFFD; (*aktu&#xFFFD; (*aktu&#xFFFD; (*aktu&#xFFFD; (*aktu&#xFFFD; (*aktu&#xFFFD; (*aktu&#xFFFD; (*aktu&#xFFFD; (*aktu&#xFFFD; (*aktu&#xFFFD; (*aktu&#xFFFD; (*aktu&#xFFFD; (*aktu&#xFFFD; (*aktu&#xFFFD; (*aktu&#xFFFD; (*aktu&#xFFFD; (*aktu&#xFFFD; (*aktu&#xFFFD; (*aktu&#xFFFD; (*aktu&#xFFFD; (*aktu&#xFFFD; (*aktu&#xFFFD; (*aktu&#xFFFD; (*aktu&#xFFFD; (*aktu&#xFFFD; (*aktu&#xFFFD; (*aktu&#xFFFD; (*aktu&#xFFFD; (*aktu&#xFFFD; (*aktu&#xFFFD; (*aktu&#xFFFD; (*aktu&#xFFFD; (*aktu&#xFFFD; (*aktu&#xFFFD; (*aktu&#xFFFD; (*aktu&#xFFFD; (*aktu&#xFFFD; (*aktu&#xFFFD; (*aktu&#xFFFD; (*aktu&#xFFFD; (*aktu&#xFFFD; (*aktu&#xFFFD; (*aktu&#xFFFD; (*aktu&#xFFFD; (*aktu&#xFFFD; (*aktu&#xFFFD; (*aktu&#xFFFD; (*aktu&#xFFFD; (*aktu&#xFFFD; (*aktu&#xFFFD; (*aktu&#xFFFD; (*aktu&#xFFFD; (*aktu&#xFFFD; (*aktu&#xFFFD; (*aktu&#xFFFD; (*aktu&#xFFFD; (*aktu&#xFFFD; (*aktu&#xFFFD; (*aktu&#xFFFD; (*aktu&#xFFFD; (*aktu&#xFFFD; (*aktu&#xFFFD; (*aktu&#xFFFD; (*aktu&#xFFFD; (*aktu&#xFFFD; (*aktu&#xFFFD; (*aktu&#xFFFD; (*aktu&#xFFFD; (*aktu&#xFFFD; (*aktu&#xFFFD; (*aktu&#xFFFD; (*aktu&#xFFFD; (*aktu&#xFFFD; (*aktu&#xFFFD; (*aktu&#xFFFD; (*aktu&#xFFFD; (*aktu&#xFFFD; (*aktu&#xFFFD; (*aktu&#xFFFD; (*aktu&#xFFFD; (*aktu&#xFFFD; (*aktu&#xFFFD; (*aktu&#xFFFD; (*aktu&#xFFFD; (*aktu&#xFFFD; (*aktu&#xFFFD; (*aktu&#xFFFD; (*aktu&#xFFFD; (*aktu&#xFFFD; (*aktu&#xFFFD; (*aktu&#xFFFD; (*aktu&#xFFFD; (*aktu&#xFFFD; (*aktu&#xFFFD; (*aktu&#xFFFD; (*aktu&#xFFFD; (*aktu&#xFFFD; (*aktu&#xFFFD; (*aktu&#xFFFD; (*aktu&#xFFFD; (*aktu&#xFFFD; (*aktu&#xFFFD; (*aktu&#xFFFD; (*aktu&#xFFFD; (*aktu&#xFFFD; (*aktu&#xFFFD; (*aktu&#xFFFD; (*aktu&#xFFFD; (*aktu&#xFFFD; (*aktu&#xFFFD; (*aktu&#xFFFD; (*aktu&#xFFFD; (*aktu&#xFFFD; (*aktu&#xFFFD; (*aktu&#xFFFD; (*aktu&#xFFFD; (*aktu&#xFFFD; (*aktu&#xFFFD; (*aktu&#xFFFD; (*aktu&#xFFFD; (*aktu&#xFFFD; (*aktu&#xFFFD; (*aktu&#xFFFD; (*aktu&#xFFFD; (*aktu&#xFFFD; (*aktu&#xFFFD; (*aktu&#xFFFD; (*aktu&#xFFFD; (*aktu&#xFFFD; (*aktu&#xFFFD; (*aktu&#xFFFD; (*aktu&#xFFFD; (*aktu&#xFFFD; (*aktu&#xFFFD; (*aktu&#xFFFD; (*aktu&#xFFFD; (*aktu&#xFFFD; (*aktu&#xFFFD; (*aktu&#xFFFD; (*aktu&#xFFFD; (*aktu&#xFFFD; (*aktu&#xFFFD; (*aktu&#xFFFD; (*aktu&#xFFFD; (*aktu&#xFFFD; (*aktu&#xFFFD; (*aktu&#xFFFD; (*aktu&#xFFFD; (*aktu&#xFFFD; (*aktu&#xFFFD; (*aktu&#xFFFD; (*aktu&#xFFFD; (*aktu&#xFFFD; (*aktu&#xFFFD; (*aktu&#xFFFD; (*aktu&#xFFFD; (*aktu&#xFFFD; (*aktu&#xFFFD; (*aktu&#xFFFD; (*aktu&#xFFFD; (*aktu&#xFFFD; (*aktu&#xFFFD; (*aktu&#xFFFD; (*aktu&#xFFFD; (*aktu&#xFFFD; (*aktu&#xFFFD; (*aktu&#xFFFD; (*aktu&#xFFFD; (*aktu&#xFFFD; (*aktu&#xFFFD; (*aktu&#xFFFD; (*aktu&#xFFFD; (*aktu&#xFFFD; (*aktu&#xFFFD; (*aktu&#xFFFD; (*aktu&#xFFFD; (*aktu&#xFFFD; (*aktu&#xFFFD; (*aktu&#xFFFD; (*aktu&#xFFFD; (*aktu&#xFFFD; (*aktu&#xFFFD; (*aktu&#xFFFD; (*aktu&#xFFFD; (*aktu&#xFFFD; (*aktu&#xFFFD; (*aktu&#xFFFD; (*aktu&#xFFFD; (*aktu&#xFFFD; (*aktu&#xFFFD; (*aktu&#xFFFD; (*aktu&#xFFFD; (*aktu&#xFFFD; (*aktu&#xFFFD; (*aktu&#xFFFD; (*aktu&#xFFFD; (*aktu&#xFFFD; (*aktu&#xFFFD; (*aktu&#xFFFD; (*aktu&#xFFFD; (*aktu&#xFFFD; (*aktu&#xFFFD; (*aktu&#xFFFD; (*aktu&#xFFFD; (*aktu&#xFFFD; (*aktu&#xFFFD; (*aktu&#xFFFD; (*aktu&#xFFFD; (*aktu&#xFFFD; (*aktu&#xFFFD; (*aktu&#xFFFD; (*aktu&#xFFFD; (*aktu&#xFFFD; (*aktu&#xFFFD; (*aktu&#xFFFD; (*aktu&#xFFFD; (*aktu&#xFFFD; (*aktu&#xFFFD; (*aktu&#xFFFD; (*aktu&#xFFFD; (*aktu&#xFFFD; (*aktu&#xFFFD; (*aktu&#xFFFD; (*aktu&#xFFFD; (*aktu&#xFFFD; (*aktu&#xFFFD; (*aktu&#xFFFD; (*aktu&#xFFFD; (*aktu&#xFFFD; (*aktu&#xFFFD; (*aktu&#xFFFD; (*aktu&#xFFFD; (*aktu&#xFFFD; (*aktu&#xFFFD; (*aktu&#xFFFD; (*aktu&#xFFFD; (*aktu&#xFFFD; (*aktu&#xFFFD; (*aktu&#xFFFD; (*aktu&#xFFFD; (*aktu&#xFFFD; (*aktu&#xFFFD; (*aktu&#xFFFD; (*aktu&#xFFFD; (*aktu&#xFFFD; (*aktu&#xFFFD; (*aktu&#xFFFD; (*aktu&#xFFFD; (*aktu&#xFFFD; (*aktu&#xFFFD; (*aktu&#xFFFD; (*aktu&#xFFFD; (*aktu&#xFFFD; (*aktu&#xFFFD; (*aktu&#xFFFD; (*aktu&#xFFFD; (*aktu&#xFFFD; (*aktu&#xFFFD; (*aktu&#xFFFD; (*aktu&#xFFFD; (*aktu&#xFFFD; (*aktu&#xFFFD; (*aktu&#xFFFD; (*aktu&#xFFFD; (*aktu&#xFFFD; (*aktu&#xFFFD; (*aktu&#xFFFD; (*aktu&#xFFFD; (*aktu&#xFFFD; (*aktu&#xFFFD; (*aktu&#xFFFD; (*aktu&#xFFFD; (*aktu&#xFFFD; (*aktu&#xFFFD; (*aktu&#xFFFD; (*aktu&#xFFFD; (*aktu&#xFFFD; (*aktu&#xFFFD; (*aktu&#xFFFD; (*aktu&#xFFFD; (*aktu&#xFFFD; (*aktu&#xFFFD; (*aktu&#xFFFD; (*aktu&#xFFFD; (*aktu&#xFFFD; (*aktu&#xFFFD; (*aktu&#xFFFD; (*aktu&#xFFFD; (*aktu&#xFFFD; (*aktu&#xFFFD; (*aktu&#xFFFD; (*aktu&#xFFFD; (*aktu&#xFFFD; (*aktu&#xFFFD; (*aktu&#xFFFD; (*aktu&#xFFFD; (*aktu&#xFFFD; (*aktu&#xFFFD; (*aktu&#xFFFD; (*aktu&#xFFFD; (*aktu&#xFFFD; (*aktu&#xFFFD; (*aktu&#xFFFD; (*aktu&#xFFFD; (*aktu&#xFFFD; (*aktu&#xFFFD; (*aktu&#xFFFD; (*aktu&#xFFFD; (*aktu&#xFFFD; (*aktu&#xFFFD; (*aktu&#xFFFD; (*aktu&#xFFFD; (*aktu&#xFFFD; (*aktu&#xFFFD; (*aktu&#xFFFD; (*aktu&#xFFFD; (*aktu&#xFFFD; (*aktu&#xFFFD; (*aktu&#xFFFD; (*aktu&#xFFFD; (*aktu&#xFFFD; (*aktu&#xFFFD; (*aktu&#xFFFD; (*aktu&#xFFFD; (*aktu&#xFFFD; (*aktu&#xFFFD; (*aktu&#xFFFD; (*aktu&#xFFFD; (*aktu&#xFFFD; (*aktu&#xFFFD; (*aktu&#xFFFD; (*aktu&#xFFFD; (*aktu&#xFFFD; (*aktu&#xFFFD; (*aktu&#xFFFD; (*aktu&#xFFFD; (*aktu&#xFFFD; (*aktu&#xFFFD; (*aktu&#xFFFD; (*aktu&#xFFFD; (*aktu&#xFFFD; (*aktu&#xFFFD; (*aktu&#xFFFD; (*aktu&#xFFFD; (*aktu&#xFFFD; (*aktu&#xFFFD; (*aktu&#xFFFD; (*aktu&#xFFFD; (*aktu&#xFFFD; (*aktu&#xFFFD; (*aktu&#xFFFD; (*aktu&#xFFFD; (*aktu&#xFFFD; (*aktu&#xFFFD; (*aktu&#xFFFD; (*aktu&#xFFFD; (*aktu&#xFFFD; (*aktu&#xFFFD; (*aktu&#xFFFD; (*aktu&#xFFFD; (*aktu&#xFFFD; (*aktu&#xFFFD; (*aktu&#xFFFD; (*aktu&#xFFFD; (*aktu&#xFFFD; (*aktu&#xFFFD; (*aktu&#xFFFD; (*aktu&#xFFFD; (*aktu&#xFFFD; (*aktu&#xFFFD; (*aktu&#xFFFD; (*aktu&#xFFFD; (*aktu&#xFFFD; (*aktu&#xFFFD; (*aktu&#xFFFD; (*aktu&#xFFFD; (*aktu&#xFFFD; (*aktu&#xFFFD; (*aktu&#xFFFD; (*aktu&#xFFFD; (*aktu&#xFFFD; (*aktu&#xFFFD; (*aktu&#xFFFD; (*aktu&#xFFFD; (*aktu&#xFFFD; (*aktu&#xFFFD; (*aktu&#xFFFD; (*aktu&#xFFFD; (*aktu&#xFFFD; (*aktu&#xFFFD; (*aktu&#xFFFD; (*aktu&#xFFFD; (*aktu&#xFFFD; (*aktu&#xFFFD; (*aktu&#xFFFD; (*aktu&#xFFFD; (*aktu&#xFFFD; (*aktu&#xFFFD; (*aktu&#xFFFD; (*aktu&#xFFFD; (*aktu&#xFFFD; (*aktu&#xFFFD; (*aktu&#xFFFD; (*aktu&#xFFFD; (*aktu&#xFFFD; (*aktu&#xFFFD; (*aktu&#xFFFD; (*aktu&#xFFFD; (*aktu&#xFFFD; (*aktu&#xFFFD; (*aktu&#xFFFD; (*aktu&#xFFFD; (*aktu&#xFFFD; (*aktu&#xFFFD; (*aktu&#xFFFD; (*aktu&#xFFFD; (*aktu&#xFFFD; (*aktu&#xFFFD; (*aktu&#xFFFD; (*aktu&#xFFFD; (*aktu&#xFFFD; (*aktu&#xFFFD; (*aktu&#xFFFD; (*aktu&#xFFFD; (*aktu&#xFFFD; (*aktu&#xFFFD; (*aktu&#xFFFD; (*aktu&#xFFFD; (*aktu&#xFFFD; (*aktu&#xFFFD; (*aktu&#xFFFD; (*aktu&#xFFFD; (*aktu&#xFFFD; (*aktu&#xFFFD; (*aktu&#xFFFD; (*aktu&#xFFFD; (*aktu&#xFFFD; (*aktu&#xFFFD; (*aktu&#xFFFD; (*aktu&#xFFFD; (*aktu&#xFFFD; (*aktu&#xFFFD; (*aktu&#xFFFD; (*aktu&#xFFFD; (*aktu&#xFFFD; (*aktu&#xFFFD; (*aktu&#xFFFD; (*aktu&#xFFFD; (*aktu&#xFFFD; (*aktu&#xFFFD; (*aktu&#xFFFD; (*aktu&#xFFFD; (*aktu&#xFFFD; (*aktu&#xFFFD; (*aktu&#xFFFD; (*aktu&#xFFFD; (*aktu&#xFFFD; (*aktu&#xFFFD; (*aktu&#xFFFD; (*aktu&#xFFFD; (*aktu&#xFFFD; (*aktu&#xFFFD; (*aktu&#xFFFD; (*aktu&#xFFFD; (*aktu&#xFFFD; (*aktu&#xFFFD; (*aktu&#xFFFD; (*aktu&#xFFFD; (*aktu&#xFFFD; (*aktu&#xFFFD; (*aktu&#xFFFD; (*aktu&#xFFFD; (*aktu&#xFFFD; (*aktu&#xFFFD; (*aktu&#xFFFD; (*aktu&#xFFFD; (*aktu&#xFFFD; (*aktu&#xFFFD; (*aktu&#xFFFD; (*aktu&#xFFFD; (*aktu&#xFFFD; (*aktu&#xFFFD; (*aktu&#xFFFD; (*aktu&#xFFFD; (*aktu&#xFFFD; (*aktu&#xFFFD; (*aktu&#xFFFD; (*aktu&#xFFFD; (*aktu&#xFFFD; (*aktu&#xFFFD; (*aktu&#xFFFD; (*aktu&#xFFFD; (*aktu&#xFFFD; (*aktu&#xFFFD; (*aktu&#xFFFD; (*aktu&#xFFFD; (*aktu&#xFFFD; (*aktu&#xFFFD; (*aktu&#xFFFD; (*aktu&#xFFFD; (*aktu&#xFFFD; (*aktu&#xFFFD; (*aktu&#xFFFD; (*aktu&#xFFFD; (*aktu&#xFFFD; (*aktu&#xFFFD; (*aktu&#xFFFD; (*aktu&#xFFFD; (*aktu&#xFFFD; (*aktu&#xFFFD; (*aktu&#xFFFD; (*aktu&#xFFFD; (*aktu&#xFFFD; (*aktu&#xFFFD; (*aktu&#xFFFD; (*aktu&#xFFFD; (*aktu&#xFFFD; (*aktu&#xFFFD; (*aktu&#xFFFD; (*aktu&#xFFFD; (*aktu&#xFFFD; (*aktu&#xFFFD; (*aktu&#xFFFD; (*aktu&#xFFFD; (*aktu&#xFFFD; (*aktu&#xFFFD; (*aktu&#xFFFD; (*aktu&#xFFFD; (*aktu&#xFFFD; (*aktu&#xFFFD; (*aktu&#xFFFD; (*aktu&#xFFFD; (*aktu&#xFFFD; (*aktu&#xFFFD; (*aktu&#xFFFD; (*aktu&#xFFFD; (*aktu&#xFFFD; (*aktu&#xFFFD; (*aktu&#xFFFD; (*aktu&#xFFFD; (*aktu&#xFFFD; (*aktu&#xFFFD; (*aktu&#xFFFD; (*aktu&#xFFFD; (*aktu&#xFFFD; (*aktu&#xFFFD; (*aktu&#xFFFD; (*aktu&#xFFFD; (*aktu&#xFFFD; (*aktu&#xFFFD; (*aktu&#xFFFD; (*aktu&#xFFFD; (*aktu&#xFFFD; (*aktu&#xFFFD; (*aktu&#xFFFD; (*aktu&#xFFFD; (*aktu&#xFFFD; (*aktu&#xFFFD; (*aktu&#xFFFD; (*aktu&#xFFFD; (*aktu&#xFFFD; (*aktu&#xFFFD; (*aktu&#xFFFD; (*aktu&#xFFFD; (*aktu&#xFFFD; (*aktu&#xFFFD; (*aktu&#xFFFD; (*aktu&#xFFFD; (*aktu&#xFFFD; (*aktu&#xFFFD; (*aktu&#xFFFD; (*aktu&#xFFFD; (*aktu&#xFFFD; (*aktu&#xFFFD; (*aktu&#xFFFD; (*aktu&#xFFFD; (*aktu&#xFFFD; (*aktu&#xFFFD; (*aktu&#xFFFD; (*aktu&#xFFFD; (*aktu&#xFFFD; (*aktu&#xFFFD; (*aktu&#xFFFD; (*aktu&#xFFFD; (*aktu&#xFFFD; (*aktu&#xFFFD; (*aktu&#xFFFD; (*aktu&#xFFFD; (*aktu&#xFFFD; (*aktu&#xFFFD; (*aktu&#xFFFD; (*aktu&#xFFFD; (*aktu&#xFFFD; (*aktu&#xFFFD; (*aktu&#xFFFD; (*aktu&#xFFFD; (*aktu&#xFFFD; (*aktu&#xFFFD; (*aktu&#xFFFD; (*aktu&#xFFFD; (*aktu&#xFFFD; (*aktu&#xFFFD; (*aktu&#xFFFD; (*aktu&#xFFFD; (*aktu&#xFFFD; (*aktu&#xFFFD; (*aktu&#xFFFD; (*aktu&#xFFFD; (*aktu&#xFFFD; (*aktu&#xFFFD; (*aktu&#xFFFD; (*aktu&#xFFFD; (*aktu&#xFFFD; (*aktu&#xFFFD; (*aktu&#xFFFD; (*aktu&#xFFFD; (*aktu&#xFFFD; (*aktu&#xFFFD; (*aktu&#xFFFD; (*aktu&#xFFFD; (*aktu&#xFFFD; (*aktu&#xFFFD; (*aktu&#xFFFD; (*aktu&#xFFFD; (*aktu&#xFFFD; (*aktu&#xFFFD; (*aktu&#xFFFD; (*aktu&#xFFFD; (*aktu&#xFFFD; (*aktu&#xFFFD;lny tlak green*)
		I_parameter :  REAL :=         0; (*parameter I PID*)
		tlak1 :  REAL :=         0; (*aktu&#xFFFD; (*aktu&#xFFFD; (*aktu&#xFFFD; (*aktu&#xFFFD; (*aktu&#xFFFD; (*aktu&#xFFFD; (*aktu&#xFFFD; (*aktu&#xFFFD; (*aktu&#xFFFD; (*aktu&#xFFFD; (*aktu&#xFFFD; (*aktu&#xFFFD; (*aktu&#xFFFD; (*aktu&#xFFFD; (*aktu&#xFFFD; (*aktu&#xFFFD; (*aktu&#xFFFD; (*aktu&#xFFFD; (*aktu&#xFFFD; (*aktu&#xFFFD; (*aktu&#xFFFD; (*aktu&#xFFFD; (*aktu&#xFFFD; (*aktu&#xFFFD; (*aktu&#xFFFD; (*aktu&#xFFFD; (*aktu&#xFFFD; (*aktu&#xFFFD; (*aktu&#xFFFD; (*aktu&#xFFFD; (*aktu&#xFFFD; (*aktu&#xFFFD; (*aktu&#xFFFD; (*aktu&#xFFFD; (*aktu&#xFFFD; (*aktu&#xFFFD; (*aktu&#xFFFD; (*aktu&#xFFFD; (*aktu&#xFFFD; (*aktu&#xFFFD; (*aktu&#xFFFD; (*aktu&#xFFFD; (*aktu&#xFFFD; (*aktu&#xFFFD; (*aktu&#xFFFD; (*aktu&#xFFFD; (*aktu&#xFFFD; (*aktu&#xFFFD; (*aktu&#xFFFD; (*aktu&#xFFFD; (*aktu&#xFFFD; (*aktu&#xFFFD; (*aktu&#xFFFD; (*aktu&#xFFFD; (*aktu&#xFFFD; (*aktu&#xFFFD; (*aktu&#xFFFD; (*aktu&#xFFFD; (*aktu&#xFFFD; (*aktu&#xFFFD; (*aktu&#xFFFD; (*aktu&#xFFFD; (*aktu&#xFFFD; (*aktu&#xFFFD; (*aktu&#xFFFD; (*aktu&#xFFFD; (*aktu&#xFFFD; (*aktu&#xFFFD; (*aktu&#xFFFD; (*aktu&#xFFFD; (*aktu&#xFFFD; (*aktu&#xFFFD; (*aktu&#xFFFD; (*aktu&#xFFFD; (*aktu&#xFFFD; (*aktu&#xFFFD; (*aktu&#xFFFD; (*aktu&#xFFFD; (*aktu&#xFFFD; (*aktu&#xFFFD; (*aktu&#xFFFD; (*aktu&#xFFFD; (*aktu&#xFFFD; (*aktu&#xFFFD; (*aktu&#xFFFD; (*aktu&#xFFFD; (*aktu&#xFFFD; (*aktu&#xFFFD; (*aktu&#xFFFD; (*aktu&#xFFFD; (*aktu&#xFFFD; (*aktu&#xFFFD; (*aktu&#xFFFD; (*aktu&#xFFFD; (*aktu&#xFFFD; (*aktu&#xFFFD; (*aktu&#xFFFD; (*aktu&#xFFFD; (*aktu&#xFFFD; (*aktu&#xFFFD; (*aktu&#xFFFD; (*aktu&#xFFFD; (*aktu&#xFFFD; (*aktu&#xFFFD; (*aktu&#xFFFD; (*aktu&#xFFFD; (*aktu&#xFFFD; (*aktu&#xFFFD; (*aktu&#xFFFD; (*aktu&#xFFFD; (*aktu&#xFFFD; (*aktu&#xFFFD; (*aktu&#xFFFD; (*aktu&#xFFFD; (*aktu&#xFFFD; (*aktu&#xFFFD; (*aktu&#xFFFD; (*aktu&#xFFFD; (*aktu&#xFFFD; (*aktu&#xFFFD; (*aktu&#xFFFD; (*aktu&#xFFFD; (*aktu&#xFFFD; (*aktu&#xFFFD; (*aktu&#xFFFD; (*aktu&#xFFFD; (*aktu&#xFFFD; (*aktu&#xFFFD; (*aktu&#xFFFD; (*aktu&#xFFFD; (*aktu&#xFFFD; (*aktu&#xFFFD; (*aktu&#xFFFD; (*aktu&#xFFFD; (*aktu&#xFFFD; (*aktu&#xFFFD; (*aktu&#xFFFD; (*aktu&#xFFFD; (*aktu&#xFFFD; (*aktu&#xFFFD; (*aktu&#xFFFD; (*aktu&#xFFFD; (*aktu&#xFFFD; (*aktu&#xFFFD; (*aktu&#xFFFD; (*aktu&#xFFFD; (*aktu&#xFFFD; (*aktu&#xFFFD; (*aktu&#xFFFD; (*aktu&#xFFFD; (*aktu&#xFFFD; (*aktu&#xFFFD; (*aktu&#xFFFD; (*aktu&#xFFFD; (*aktu&#xFFFD; (*aktu&#xFFFD; (*aktu&#xFFFD; (*aktu&#xFFFD; (*aktu&#xFFFD; (*aktu&#xFFFD; (*aktu&#xFFFD; (*aktu&#xFFFD; (*aktu&#xFFFD; (*aktu&#xFFFD; (*aktu&#xFFFD; (*aktu&#xFFFD; (*aktu&#xFFFD; (*aktu&#xFFFD; (*aktu&#xFFFD; (*aktu&#xFFFD; (*aktu&#xFFFD; (*aktu&#xFFFD; (*aktu&#xFFFD; (*aktu&#xFFFD; (*aktu&#xFFFD; (*aktu&#xFFFD; (*aktu&#xFFFD; (*aktu&#xFFFD; (*aktu&#xFFFD; (*aktu&#xFFFD; (*aktu&#xFFFD; (*aktu&#xFFFD; (*aktu&#xFFFD; (*aktu&#xFFFD; (*aktu&#xFFFD; (*aktu&#xFFFD; (*aktu&#xFFFD; (*aktu&#xFFFD; (*aktu&#xFFFD; (*aktu&#xFFFD; (*aktu&#xFFFD; (*aktu&#xFFFD; (*aktu&#xFFFD; (*aktu&#xFFFD; (*aktu&#xFFFD; (*aktu&#xFFFD; (*aktu&#xFFFD; (*aktu&#xFFFD; (*aktu&#xFFFD; (*aktu&#xFFFD; (*aktu&#xFFFD; (*aktu&#xFFFD; (*aktu&#xFFFD; (*aktu&#xFFFD; (*aktu&#xFFFD; (*aktu&#xFFFD; (*aktu&#xFFFD; (*aktu&#xFFFD; (*aktu&#xFFFD; (*aktu&#xFFFD; (*aktu&#xFFFD; (*aktu&#xFFFD; (*aktu&#xFFFD; (*aktu&#xFFFD; (*aktu&#xFFFD; (*aktu&#xFFFD; (*aktu&#xFFFD; (*aktu&#xFFFD; (*aktu&#xFFFD; (*aktu&#xFFFD; (*aktu&#xFFFD; (*aktu&#xFFFD; (*aktu&#xFFFD; (*aktu&#xFFFD; (*aktu&#xFFFD; (*aktu&#xFFFD; (*aktu&#xFFFD; (*aktu&#xFFFD; (*aktu&#xFFFD; (*aktu&#xFFFD; (*aktu&#xFFFD; (*aktu&#xFFFD; (*aktu&#xFFFD; (*aktu&#xFFFD; (*aktu&#xFFFD; (*aktu&#xFFFD; (*aktu&#xFFFD; (*aktu&#xFFFD; (*aktu&#xFFFD; (*aktu&#xFFFD; (*aktu&#xFFFD; (*aktu&#xFFFD; (*aktu&#xFFFD; (*aktu&#xFFFD; (*aktu&#xFFFD; (*aktu&#xFFFD; (*aktu&#xFFFD; (*aktu&#xFFFD; (*aktu&#xFFFD; (*aktu&#xFFFD; (*aktu&#xFFFD; (*aktu&#xFFFD; (*aktu&#xFFFD; (*aktu&#xFFFD; (*aktu&#xFFFD; (*aktu&#xFFFD; (*aktu&#xFFFD; (*aktu&#xFFFD; (*aktu&#xFFFD; (*aktu&#xFFFD; (*aktu&#xFFFD; (*aktu&#xFFFD; (*aktu&#xFFFD; (*aktu&#xFFFD; (*aktu&#xFFFD; (*aktu&#xFFFD; (*aktu&#xFFFD; (*aktu&#xFFFD; (*aktu&#xFFFD; (*aktu&#xFFFD; (*aktu&#xFFFD; (*aktu&#xFFFD; (*aktu&#xFFFD; (*aktu&#xFFFD; (*aktu&#xFFFD; (*aktu&#xFFFD; (*aktu&#xFFFD; (*aktu&#xFFFD; (*aktu&#xFFFD; (*aktu&#xFFFD; (*aktu&#xFFFD; (*aktu&#xFFFD; (*aktu&#xFFFD; (*aktu&#xFFFD; (*aktu&#xFFFD; (*aktu&#xFFFD; (*aktu&#xFFFD; (*aktu&#xFFFD; (*aktu&#xFFFD; (*aktu&#xFFFD; (*aktu&#xFFFD; (*aktu&#xFFFD; (*aktu&#xFFFD; (*aktu&#xFFFD; (*aktu&#xFFFD; (*aktu&#xFFFD; (*aktu&#xFFFD; (*aktu&#xFFFD; (*aktu&#xFFFD; (*aktu&#xFFFD; (*aktu&#xFFFD; (*aktu&#xFFFD; (*aktu&#xFFFD; (*aktu&#xFFFD; (*aktu&#xFFFD; (*aktu&#xFFFD; (*aktu&#xFFFD; (*aktu&#xFFFD; (*aktu&#xFFFD; (*aktu&#xFFFD; (*aktu&#xFFFD; (*aktu&#xFFFD; (*aktu&#xFFFD; (*aktu&#xFFFD; (*aktu&#xFFFD; (*aktu&#xFFFD; (*aktu&#xFFFD; (*aktu&#xFFFD; (*aktu&#xFFFD; (*aktu&#xFFFD; (*aktu&#xFFFD; (*aktu&#xFFFD; (*aktu&#xFFFD; (*aktu&#xFFFD; (*aktu&#xFFFD; (*aktu&#xFFFD; (*aktu&#xFFFD; (*aktu&#xFFFD; (*aktu&#xFFFD; (*aktu&#xFFFD; (*aktu&#xFFFD; (*aktu&#xFFFD; (*aktu&#xFFFD; (*aktu&#xFFFD; (*aktu&#xFFFD; (*aktu&#xFFFD; (*aktu&#xFFFD; (*aktu&#xFFFD; (*aktu&#xFFFD; (*aktu&#xFFFD; (*aktu&#xFFFD; (*aktu&#xFFFD; (*aktu&#xFFFD; (*aktu&#xFFFD; (*aktu&#xFFFD; (*aktu&#xFFFD; (*aktu&#xFFFD; (*aktu&#xFFFD; (*aktu&#xFFFD; (*aktu&#xFFFD; (*aktu&#xFFFD; (*aktu&#xFFFD; (*aktu&#xFFFD; (*aktu&#xFFFD; (*aktu&#xFFFD; (*aktu&#xFFFD; (*aktu&#xFFFD; (*aktu&#xFFFD; (*aktu&#xFFFD; (*aktu&#xFFFD; (*aktu&#xFFFD; (*aktu&#xFFFD; (*aktu&#xFFFD; (*aktu&#xFFFD; (*aktu&#xFFFD; (*aktu&#xFFFD; (*aktu&#xFFFD; (*aktu&#xFFFD; (*aktu&#xFFFD; (*aktu&#xFFFD; (*aktu&#xFFFD; (*aktu&#xFFFD; (*aktu&#xFFFD; (*aktu&#xFFFD; (*aktu&#xFFFD; (*aktu&#xFFFD; (*aktu&#xFFFD; (*aktu&#xFFFD; (*aktu&#xFFFD; (*aktu&#xFFFD; (*aktu&#xFFFD; (*aktu&#xFFFD; (*aktu&#xFFFD; (*aktu&#xFFFD; (*aktu&#xFFFD; (*aktu&#xFFFD; (*aktu&#xFFFD; (*aktu&#xFFFD; (*aktu&#xFFFD; (*aktu&#xFFFD; (*aktu&#xFFFD; (*aktu&#xFFFD; (*aktu&#xFFFD; (*aktu&#xFFFD; (*aktu&#xFFFD; (*aktu&#xFFFD; (*aktu&#xFFFD; (*aktu&#xFFFD; (*aktu&#xFFFD; (*aktu&#xFFFD; (*aktu&#xFFFD; (*aktu&#xFFFD; (*aktu&#xFFFD; (*aktu&#xFFFD; (*aktu&#xFFFD; (*aktu&#xFFFD; (*aktu&#xFFFD; (*aktu&#xFFFD; (*aktu&#xFFFD; (*aktu&#xFFFD; (*aktu&#xFFFD; (*aktu&#xFFFD; (*aktu&#xFFFD; (*aktu&#xFFFD; (*aktu&#xFFFD; (*aktu&#xFFFD; (*aktu&#xFFFD; (*aktu&#xFFFD; (*aktu&#xFFFD; (*aktu&#xFFFD; (*aktu&#xFFFD; (*aktu&#xFFFD; (*aktu&#xFFFD; (*aktu&#xFFFD; (*aktu&#xFFFD; (*aktu&#xFFFD; (*aktu&#xFFFD; (*aktu&#xFFFD; (*aktu&#xFFFD; (*aktu&#xFFFD; (*aktu&#xFFFD; (*aktu&#xFFFD; (*aktu&#xFFFD; (*aktu&#xFFFD; (*aktu&#xFFFD; (*aktu&#xFFFD; (*aktu&#xFFFD; (*aktu&#xFFFD; (*aktu&#xFFFD; (*aktu&#xFFFD; (*aktu&#xFFFD; (*aktu&#xFFFD; (*aktu&#xFFFD; (*aktu&#xFFFD; (*aktu&#xFFFD; (*aktu&#xFFFD; (*aktu&#xFFFD; (*aktu&#xFFFD; (*aktu&#xFFFD; (*aktu&#xFFFD; (*aktu&#xFFFD; (*aktu&#xFFFD; (*aktu&#xFFFD; (*aktu&#xFFFD; (*aktu&#xFFFD; (*aktu&#xFFFD; (*aktu&#xFFFD; (*aktu&#xFFFD; (*aktu&#xFFFD; (*aktu&#xFFFD; (*aktu&#xFFFD; (*aktu&#xFFFD; (*aktu&#xFFFD; (*aktu&#xFFFD; (*aktu&#xFFFD; (*aktu&#xFFFD; (*aktu&#xFFFD; (*aktu&#xFFFD; (*aktu&#xFFFD; (*aktu&#xFFFD; (*aktu&#xFFFD; (*aktu&#xFFFD; (*aktu&#xFFFD; (*aktu&#xFFFD; (*aktu&#xFFFD; (*aktu&#xFFFD; (*aktu&#xFFFD; (*aktu&#xFFFD; (*aktu&#xFFFD; (*aktu&#xFFFD; (*aktu&#xFFFD; (*aktu&#xFFFD; (*aktu&#xFFFD; (*aktu&#xFFFD; (*aktu&#xFFFD; (*aktu&#xFFFD; (*aktu&#xFFFD; (*aktu&#xFFFD; (*aktu&#xFFFD; (*aktu&#xFFFD; (*aktu&#xFFFD; (*aktu&#xFFFD; (*aktu&#xFFFD; (*aktu&#xFFFD; (*aktu&#xFFFD; (*aktu&#xFFFD; (*aktu&#xFFFD; (*aktu&#xFFFD; (*aktu&#xFFFD; (*aktu&#xFFFD; (*aktu&#xFFFD; (*aktu&#xFFFD; (*aktu&#xFFFD; (*aktu&#xFFFD; (*aktu&#xFFFD; (*aktu&#xFFFD; (*aktu&#xFFFD; (*aktu&#xFFFD; (*aktu&#xFFFD; (*aktu&#xFFFD; (*aktu&#xFFFD; (*aktu&#xFFFD; (*aktu&#xFFFD; (*aktu&#xFFFD; (*aktu&#xFFFD; (*aktu&#xFFFD; (*aktu&#xFFFD; (*aktu&#xFFFD; (*aktu&#xFFFD; (*aktu&#xFFFD; (*aktu&#xFFFD; (*aktu&#xFFFD; (*aktu&#xFFFD; (*aktu&#xFFFD; (*aktu&#xFFFD; (*aktu&#xFFFD; (*aktu&#xFFFD; (*aktu&#xFFFD; (*aktu&#xFFFD; (*aktu&#xFFFD; (*aktu&#xFFFD; (*aktu&#xFFFD; (*aktu&#xFFFD; (*aktu&#xFFFD; (*aktu&#xFFFD; (*aktu&#xFFFD; (*aktu&#xFFFD; (*aktu&#xFFFD; (*aktu&#xFFFD; (*aktu&#xFFFD; (*aktu&#xFFFD; (*aktu&#xFFFD; (*aktu&#xFFFD; (*aktu&#xFFFD; (*aktu&#xFFFD; (*aktu&#xFFFD; (*aktu&#xFFFD; (*aktu&#xFFFD; (*aktu&#xFFFD; (*aktu&#xFFFD; (*aktu&#xFFFD; (*aktu&#xFFFD; (*aktu&#xFFFD; (*aktu&#xFFFD; (*aktu&#xFFFD; (*aktu&#xFFFD; (*aktu&#xFFFD; (*aktu&#xFFFD; (*aktu&#xFFFD; (*aktu&#xFFFD; (*aktu&#xFFFD; (*aktu&#xFFFD; (*aktu&#xFFFD; (*aktu&#xFFFD; (*aktu&#xFFFD; (*aktu&#xFFFD; (*aktu&#xFFFD; (*aktu&#xFFFD; (*aktu&#xFFFD; (*aktu&#xFFFD; (*aktu&#xFFFD; (*aktu&#xFFFD; (*aktu&#xFFFD; (*aktu&#xFFFD; (*aktu&#xFFFD; (*aktu&#xFFFD; (*aktu&#xFFFD; (*aktu&#xFFFD; (*aktu&#xFFFD; (*aktu&#xFFFD; (*aktu&#xFFFD; (*aktu&#xFFFD; (*aktu&#xFFFD; (*aktu&#xFFFD; (*aktu&#xFFFD; (*aktu&#xFFFD; (*aktu&#xFFFD; (*aktu&#xFFFD; (*aktu&#xFFFD; (*aktu&#xFFFD; (*aktu&#xFFFD; (*aktu&#xFFFD; (*aktu&#xFFFD; (*aktu&#xFFFD; (*aktu&#xFFFD; (*aktu&#xFFFD; (*aktu&#xFFFD; (*aktu&#xFFFD; (*aktu&#xFFFD; (*aktu&#xFFFD; (*aktu&#xFFFD; (*aktu&#xFFFD; (*aktu&#xFFFD; (*aktu&#xFFFD; (*aktu&#xFFFD; (*aktu&#xFFFD; (*aktu&#xFFFD; (*aktu&#xFFFD; (*aktu&#xFFFD; (*aktu&#xFFFD; (*aktu&#xFFFD; (*aktu&#xFFFD; (*aktu&#xFFFD; (*aktu&#xFFFD; (*aktu&#xFFFD; (*aktu&#xFFFD; (*aktu&#xFFFD; (*aktu&#xFFFD; (*aktu&#xFFFD; (*aktu&#xFFFD; (*aktu&#xFFFD; (*aktu&#xFFFD; (*aktu&#xFFFD; (*aktu&#xFFFD; (*aktu&#xFFFD; (*aktu&#xFFFD; (*aktu&#xFFFD; (*aktu&#xFFFD; (*aktu&#xFFFD; (*aktu&#xFFFD; (*aktu&#xFFFD; (*aktu&#xFFFD; (*aktu&#xFFFD; (*aktu&#xFFFD; (*aktu&#xFFFD; (*aktu&#xFFFD; (*aktu&#xFFFD; (*aktu&#xFFFD; (*aktu&#xFFFD; (*aktu&#xFFFD; (*aktu&#xFFFD; (*aktu&#xFFFD; (*aktu&#xFFFD; (*aktu&#xFFFD; (*aktu&#xFFFD; (*aktu&#xFFFD; (*aktu&#xFFFD; (*aktu&#xFFFD; (*aktu&#xFFFD; (*aktu&#xFFFD; (*aktu&#xFFFD; (*aktu&#xFFFD; (*aktu&#xFFFD; (*aktu&#xFFFD; (*aktu&#xFFFD; (*aktu&#xFFFD; (*aktu&#xFFFD; (*aktu&#xFFFD; (*aktu&#xFFFD; (*aktu&#xFFFD; (*aktu&#xFFFD; (*aktu&#xFFFD; (*aktu&#xFFFD; (*aktu&#xFFFD; (*aktu&#xFFFD; (*aktu&#xFFFD; (*aktu&#xFFFD; (*aktu&#xFFFD; (*aktu&#xFFFD; (*aktu&#xFFFD; (*aktu&#xFFFD; (*aktu&#xFFFD; (*aktu&#xFFFD; (*aktu&#xFFFD; (*aktu&#xFFFD; (*aktu&#xFFFD; (*aktu&#xFFFD; (*aktu&#xFFFD; (*aktu&#xFFFD; (*aktu&#xFFFD; (*aktu&#xFFFD; (*aktu&#xFFFD; (*aktu&#xFFFD; (*aktu&#xFFFD; (*aktu&#xFFFD; (*aktu&#xFFFD; (*aktu&#xFFFD; (*aktu&#xFFFD; (*aktu&#xFFFD; (*aktu&#xFFFD; (*aktu&#xFFFD; (*aktu&#xFFFD; (*aktu&#xFFFD; (*aktu&#xFFFD; (*aktu&#xFFFD; (*aktu&#xFFFD; (*aktu&#xFFFD; (*aktu&#xFFFD; (*aktu&#xFFFD; (*aktu&#xFFFD; (*aktu&#xFFFD; (*aktu&#xFFFD; (*aktu&#xFFFD; (*aktu&#xFFFD; (*aktu&#xFFFD; (*aktu&#xFFFD; (*aktu&#xFFFD; (*aktu&#xFFFD; (*aktu&#xFFFD; (*aktu&#xFFFD; (*aktu&#xFFFD; (*aktu&#xFFFD; (*aktu&#xFFFD; (*aktu&#xFFFD; (*aktu&#xFFFD; (*aktu&#xFFFD; (*aktu&#xFFFD; (*aktu&#xFFFD; (*aktu&#xFFFD; (*aktu&#xFFFD; (*aktu&#xFFFD; (*aktu&#xFFFD; (*aktu&#xFFFD; (*aktu&#xFFFD; (*aktu&#xFFFD; (*aktu&#xFFFD; (*aktu&#xFFFD; (*aktu&#xFFFD; (*aktu&#xFFFD; (*aktu&#xFFFD; (*aktu&#xFFFD; (*aktu&#xFFFD; (*aktu&#xFFFD; (*aktu&#xFFFD; (*aktu&#xFFFD; (*aktu&#xFFFD; (*aktu&#xFFFD; (*aktu&#xFFFD; (*aktu&#xFFFD; (*aktu&#xFFFD; (*aktu&#xFFFD; (*aktu&#xFFFD; (*aktu&#xFFFD; (*aktu&#xFFFD; (*aktu&#xFFFD; (*aktu&#xFFFD; (*aktu&#xFFFD; (*aktu&#xFFFD; (*aktu&#xFFFD; (*aktu&#xFFFD; (*aktu&#xFFFD; (*aktu&#xFFFD; (*aktu&#xFFFD; (*aktu&#xFFFD; (*aktu&#xFFFD; (*aktu&#xFFFD; (*aktu&#xFFFD; (*aktu&#xFFFD; (*aktu&#xFFFD; (*aktu&#xFFFD; (*aktu&#xFFFD; (*aktu&#xFFFD; (*aktu&#xFFFD; (*aktu&#xFFFD; (*aktu&#xFFFD; (*aktu&#xFFFD; (*aktu&#xFFFD; (*aktu&#xFFFD; (*aktu&#xFFFD; (*aktu&#xFFFD; (*aktu&#xFFFD; (*aktu&#xFFFD; (*aktu&#xFFFD; (*aktu&#xFFFD; (*aktu&#xFFFD; (*aktu&#xFFFD; (*aktu&#xFFFD; (*aktu&#xFFFD; (*aktu&#xFFFD; (*aktu&#xFFFD; (*aktu&#xFFFD; (*aktu&#xFFFD; (*aktu&#xFFFD; (*aktu&#xFFFD; (*aktu&#xFFFD; (*aktu&#xFFFD; (*aktu&#xFFFD; (*aktu&#xFFFD; (*aktu&#xFFFD; (*aktu&#xFFFD; (*aktu&#xFFFD; (*aktu&#xFFFD; (*aktu&#xFFFD; (*aktu&#xFFFD; (*aktu&#xFFFD; (*aktu&#xFFFD; (*aktu&#xFFFD; (*aktu&#xFFFD; (*aktu&#xFFFD; (*aktu&#xFFFD; (*aktu&#xFFFD; (*aktu&#xFFFD; (*aktu&#xFFFD; (*aktu&#xFFFD; (*aktu&#xFFFD; (*aktu&#xFFFD; (*aktu&#xFFFD; (*aktu&#xFFFD; (*aktu&#xFFFD; (*aktu&#xFFFD; (*aktu&#xFFFD; (*aktu&#xFFFD; (*aktu&#xFFFD; (*aktu&#xFFFD; (*aktu&#xFFFD; (*aktu&#xFFFD; (*aktu&#xFFFD; (*aktu&#xFFFD; (*aktu&#xFFFD; (*aktu&#xFFFD; (*aktu&#xFFFD; (*aktu&#xFFFD; (*aktu&#xFFFD; (*aktu&#xFFFD; (*aktu&#xFFFD; (*aktu&#xFFFD; (*aktu&#xFFFD; (*aktu&#xFFFD; (*aktu&#xFFFD; (*aktu&#xFFFD; (*aktu&#xFFFD; (*aktu&#xFFFD; (*aktu&#xFFFD; (*aktu&#xFFFD; (*aktu&#xFFFD; (*aktu&#xFFFD; (*aktu&#xFFFD; (*aktu&#xFFFD; (*aktu&#xFFFD; (*aktu&#xFFFD; (*aktu&#xFFFD; (*aktu&#xFFFD; (*aktu&#xFFFD; (*aktu&#xFFFD; (*aktu&#xFFFD; (*aktu&#xFFFD; (*aktu&#xFFFD; (*aktu&#xFFFD; (*aktu&#xFFFD; (*aktu&#xFFFD; (*aktu&#xFFFD; (*aktu&#xFFFD; (*aktu&#xFFFD; (*aktu&#xFFFD; (*aktu&#xFFFD; (*aktu&#xFFFD; (*aktu&#xFFFD; (*aktu&#xFFFD; (*aktu&#xFFFD; (*aktu&#xFFFD; (*aktu&#xFFFD; (*aktu&#xFFFD; (*aktu&#xFFFD; (*aktu&#xFFFD; (*aktu&#xFFFD; (*aktu&#xFFFD; (*aktu&#xFFFD; (*aktu&#xFFFD; (*aktu&#xFFFD; (*aktu&#xFFFD; (*aktu&#xFFFD; (*aktu&#xFFFD; (*aktu&#xFFFD; (*aktu&#xFFFD; (*aktu&#xFFFD; (*aktu&#xFFFD; (*aktu&#xFFFD; (*aktu&#xFFFD; (*aktu&#xFFFD; (*aktu&#xFFFD; (*aktu&#xFFFD; (*aktu&#xFFFD; (*aktu&#xFFFD; (*aktu&#xFFFD; (*aktu&#xFFFD; (*aktu&#xFFFD; (*aktu&#xFFFD; (*aktu&#xFFFD; (*aktu&#xFFFD; (*aktu&#xFFFD; (*aktu&#xFFFD; (*aktu&#xFFFD; (*aktu&#xFFFD; (*aktu&#xFFFD; (*aktu&#xFFFD; (*aktu&#xFFFD; (*aktu&#xFFFD; (*aktu&#xFFFD; (*aktu&#xFFFD; (*aktu&#xFFFD; (*aktu&#xFFFD; (*aktu&#xFFFD; (*aktu&#xFFFD; (*aktu&#xFFFD; (*aktu&#xFFFD; (*aktu&#xFFFD; (*aktu&#xFFFD; (*aktu&#xFFFD; (*aktu&#xFFFD; (*aktu&#xFFFD; (*aktu&#xFFFD; (*aktu&#xFFFD; (*aktu&#xFFFD; (*aktu&#xFFFD; (*aktu&#xFFFD; (*aktu&#xFFFD; (*aktu&#xFFFD; (*aktu&#xFFFD; (*aktu&#xFFFD; (*aktu&#xFFFD; (*aktu&#xFFFD; (*aktu&#xFFFD; (*aktu&#xFFFD; (*aktu&#xFFFD; (*aktu&#xFFFD; (*aktu&#xFFFD; (*aktu&#xFFFD; (*aktu&#xFFFD; (*aktu&#xFFFD; (*aktu&#xFFFD; (*aktu&#xFFFD; (*aktu&#xFFFD; (*aktu&#xFFFD; (*aktu&#xFFFD; (*aktu&#xFFFD; (*aktu&#xFFFD; (*aktu&#xFFFD; (*aktu&#xFFFD; (*aktu&#xFFFD; (*aktu&#xFFFD; (*aktu&#xFFFD; (*aktu&#xFFFD; (*aktu&#xFFFD; (*aktu&#xFFFD; (*aktu&#xFFFD; (*aktu&#xFFFD; (*aktu&#xFFFD; (*aktu&#xFFFD; (*aktu&#xFFFD; (*aktu&#xFFFD; (*aktu&#xFFFD; (*aktu&#xFFFD; (*aktu&#xFFFD; (*aktu&#xFFFD; (*aktu&#xFFFD; (*aktu&#xFFFD; (*aktu&#xFFFD; (*aktu&#xFFFD; (*aktu&#xFFFD; (*aktu&#xFFFD; (*aktu&#xFFFD; (*aktu&#xFFFD; (*aktu&#xFFFD; (*aktu&#xFFFD; (*aktu&#xFFFD; (*aktu&#xFFFD; (*aktu&#xFFFD; (*aktu&#xFFFD; (*aktu&#xFFFD; (*aktu&#xFFFD; (*aktu&#xFFFD; (*aktu&#xFFFD; (*aktu&#xFFFD; (*aktu&#xFFFD; (*aktu&#xFFFD; (*aktu&#xFFFD; (*aktu&#xFFFD; (*aktu&#xFFFD; (*aktu&#xFFFD; (*aktu&#xFFFD; (*aktu&#xFFFD; (*aktu&#xFFFD; (*aktu&#xFFFD; (*aktu&#xFFFD; (*aktu&#xFFFD; (*aktu&#xFFFD; (*aktu&#xFFFD; (*aktu&#xFFFD; (*aktu&#xFFFD; (*aktu&#xFFFD; (*aktu&#xFFFD; (*aktu&#xFFFD; (*aktu&#xFFFD; (*aktu&#xFFFD; (*aktu&#xFFFD; (*aktu&#xFFFD; (*aktu&#xFFFD; (*aktu&#xFFFD; (*aktu&#xFFFD; (*aktu&#xFFFD; (*aktu&#xFFFD; (*aktu&#xFFFD; (*aktu&#xFFFD; (*aktu&#xFFFD; (*aktu&#xFFFD; (*aktu&#xFFFD; (*aktu&#xFFFD; (*aktu&#xFFFD; (*aktu&#xFFFD; (*aktu&#xFFFD; (*aktu&#xFFFD; (*aktu&#xFFFD; (*aktu&#xFFFD; (*aktu&#xFFFD; (*aktu&#xFFFD; (*aktu&#xFFFD; (*aktu&#xFFFD; (*aktu&#xFFFD; (*aktu&#xFFFD; (*aktu&#xFFFD; (*aktu&#xFFFD; (*aktu&#xFFFD; (*aktu&#xFFFD; (*aktu&#xFFFD; (*aktu&#xFFFD; (*aktu&#xFFFD; (*aktu&#xFFFD; (*aktu&#xFFFD; (*aktu&#xFFFD; (*aktu&#xFFFD; (*aktu&#xFFFD; (*aktu&#xFFFD; (*aktu&#xFFFD; (*aktu&#xFFFD; (*aktu&#xFFFD; (*aktu&#xFFFD; (*aktu&#xFFFD; (*aktu&#xFFFD; (*aktu&#xFFFD; (*aktu&#xFFFD; (*aktu&#xFFFD; (*aktu&#xFFFD; (*aktu&#xFFFD; (*aktu&#xFFFD; (*aktu&#xFFFD; (*aktu&#xFFFD; (*aktu&#xFFFD; (*aktu&#xFFFD; (*aktu&#xFFFD; (*aktu&#xFFFD; (*aktu&#xFFFD; (*aktu&#xFFFD; (*aktu&#xFFFD; (*aktu&#xFFFD; (*aktu&#xFFFD; (*aktu&#xFFFD; (*aktu&#xFFFD; (*aktu&#xFFFD; (*aktu&#xFFFD; (*aktu&#xFFFD; (*aktu&#xFFFD; (*aktu&#xFFFD; (*aktu&#xFFFD; (*aktu&#xFFFD; (*aktu&#xFFFD; (*aktu&#xFFFD; (*aktu&#xFFFD; (*aktu&#xFFFD; (*aktu&#xFFFD; (*aktu&#xFFFD; (*aktu&#xFFFD; (*aktu&#xFFFD; (*aktu&#xFFFD; (*aktu&#xFFFD; (*aktu&#xFFFD; (*aktu&#xFFFD; (*aktu&#xFFFD; (*aktu&#xFFFD; (*aktu&#xFFFD; (*aktu&#xFFFD; (*aktu&#xFFFD; (*aktu&#xFFFD; (*aktu&#xFFFD; (*aktu&#xFFFD; (*aktu&#xFFFD; (*aktu&#xFFFD; (*aktu&#xFFFD; (*aktu&#xFFFD; (*aktu&#xFFFD; (*aktu&#xFFFD; (*aktu&#xFFFD; (*aktu&#xFFFD; (*aktu&#xFFFD; (*aktu&#xFFFD; (*aktu&#xFFFD; (*aktu&#xFFFD; (*aktu&#xFFFD; (*aktu&#xFFFD; (*aktu&#xFFFD; (*aktu&#xFFFD; (*aktu&#xFFFD; (*aktu&#xFFFD; (*aktu&#xFFFD; (*aktu&#xFFFD; (*aktu&#xFFFD; (*aktu&#xFFFD; (*aktu&#xFFFD; (*aktu&#xFFFD; (*aktu&#xFFFD; (*aktu&#xFFFD; (*aktu&#xFFFD; (*aktu&#xFFFD; (*aktu&#xFFFD; (*aktu&#xFFFD; (*aktu&#xFFFD; (*aktu&#xFFFD; (*aktu&#xFFFD; (*aktu&#xFFFD; (*aktu&#xFFFD; (*aktu&#xFFFD; (*aktu&#xFFFD; (*aktu&#xFFFD; (*aktu&#xFFFD; (*aktu&#xFFFD; (*aktu&#xFFFD; (*aktu&#xFFFD; (*aktu&#xFFFD; (*aktu&#xFFFD; (*aktu&#xFFFD; (*aktu&#xFFFD; (*aktu&#xFFFD; (*aktu&#xFFFD; (*aktu&#xFFFD; (*aktu&#xFFFD; (*aktu&#xFFFD; (*aktu&#xFFFD; (*aktu&#xFFFD; (*aktu&#xFFFD; (*aktu&#xFFFD; (*aktu&#xFFFD; (*aktu&#xFFFD; (*aktu&#xFFFD; (*aktu&#xFFFD; (*aktu&#xFFFD; (*aktu&#xFFFD; (*aktu&#xFFFD; (*aktu&#xFFFD; (*aktu&#xFFFD; (*aktu&#xFFFD; (*aktu&#xFFFD; (*aktu&#xFFFD; (*aktu&#xFFFD; (*aktu&#xFFFD; (*aktu&#xFFFD; (*aktu&#xFFFD; (*aktu&#xFFFD; (*aktu&#xFFFD; (*aktu&#xFFFD; (*aktu&#xFFFD; (*aktu&#xFFFD; (*aktu&#xFFFD; (*aktu&#xFFFD; (*aktu&#xFFFD; (*aktu&#xFFFD; (*aktu&#xFFFD; (*aktu&#xFFFD; (*aktu&#xFFFD; (*aktu&#xFFFD; (*aktu&#xFFFD; (*aktu&#xFFFD; (*aktu&#xFFFD; (*aktu&#xFFFD; (*aktu&#xFFFD; (*aktu&#xFFFD; (*aktu&#xFFFD; (*aktu&#xFFFD; (*aktu&#xFFFD; (*aktu&#xFFFD; (*aktu&#xFFFD; (*aktu&#xFFFD; (*aktu&#xFFFD; (*aktu&#xFFFD; (*aktu&#xFFFD; (*aktu&#xFFFD; (*aktu&#xFFFD; (*aktu&#xFFFD; (*aktu&#xFFFD; (*aktu&#xFFFD; (*aktu&#xFFFD; (*aktu&#xFFFD; (*aktu&#xFFFD; (*aktu&#xFFFD; (*aktu&#xFFFD; (*aktu&#xFFFD; (*aktu&#xFFFD; (*aktu&#xFFFD; (*aktu&#xFFFD; (*aktu&#xFFFD; (*aktu&#xFFFD; (*aktu&#xFFFD; (*aktu&#xFFFD; (*aktu&#xFFFD; (*aktu&#xFFFD; (*aktu&#xFFFD; (*aktu&#xFFFD; (*aktu&#xFFFD; (*aktu&#xFFFD; (*aktu&#xFFFD; (*aktu&#xFFFD; (*aktu&#xFFFD; (*aktu&#xFFFD; (*aktu&#xFFFD; (*aktu&#xFFFD; (*aktu&#xFFFD; (*aktu&#xFFFD; (*aktu&#xFFFD; (*aktu&#xFFFD; (*aktu&#xFFFD; (*aktu&#xFFFD; (*aktu&#xFFFD; (*aktu&#xFFFD; (*aktu&#xFFFD; (*aktu&#xFFFD; (*aktu&#xFFFD; (*aktu&#xFFFD; (*aktu&#xFFFD; (*aktu&#xFFFD; (*aktu&#xFFFD; (*aktu&#xFFFD; (*aktu&#xFFFD; (*aktu&#xFFFD; (*aktu&#xFFFD; (*aktu&#xFFFD; (*aktu&#xFFFD; (*aktu&#xFFFD; (*aktu&#xFFFD; (*aktu&#xFFFD; (*aktu&#xFFFD; (*aktu&#xFFFD; (*aktu&#xFFFD; (*aktu&#xFFFD; (*aktu&#xFFFD; (*aktu&#xFFFD; (*aktu&#xFFFD; (*aktu&#xFFFD; (*aktu&#xFFFD; (*aktu&#xFFFD; (*aktu&#xFFFD; (*aktu&#xFFFD; (*aktu&#xFFFD; (*aktu&#xFFFD; (*aktu&#xFFFD; (*aktu&#xFFFD; (*aktu&#xFFFD; (*aktu&#xFFFD; (*aktu&#xFFFD; (*aktu&#xFFFD; (*aktu&#xFFFD; (*aktu&#xFFFD; (*aktu&#xFFFD; (*aktu&#xFFFD; (*aktu&#xFFFD; (*aktu&#xFFFD; (*aktu&#xFFFD; (*aktu&#xFFFD; (*aktu&#xFFFD; (*aktu&#xFFFD; (*aktu&#xFFFD; (*aktu&#xFFFD; (*aktu&#xFFFD; (*aktu&#xFFFD; (*aktu&#xFFFD; (*aktu&#xFFFD; (*aktu&#xFFFD; (*aktu&#xFFFD; (*aktu&#xFFFD; (*aktu&#xFFFD; (*aktu&#xFFFD; (*aktu&#xFFFD; (*aktu&#xFFFD; (*aktu&#xFFFD; (*aktu&#xFFFD; (*aktu&#xFFFD; (*aktu&#xFFFD; (*aktu&#xFFFD; (*aktu&#xFFFD; (*aktu&#xFFFD; (*aktu&#xFFFD; (*aktu&#xFFFD; (*aktu&#xFFFD; (*aktu&#xFFFD; (*aktu&#xFFFD; (*aktu&#xFFFD; (*aktu&#xFFFD; (*aktu&#xFFFD; (*aktu&#xFFFD; (*aktu&#xFFFD; (*aktu&#xFFFD; (*aktu&#xFFFD; (*aktu&#xFFFD; (*aktu&#xFFFD; (*aktu&#xFFFD; (*aktu&#xFFFD; (*aktu&#xFFFD; (*aktu&#xFFFD; (*aktu&#xFFFD; (*aktu&#xFFFD; (*aktu&#xFFFD; (*aktu&#xFFFD; (*aktu&#xFFFD; (*aktu&#xFFFD; (*aktu&#xFFFD; (*aktu&#xFFFD; (*aktu&#xFFFD; (*aktu&#xFFFD; (*aktu&#xFFFD; (*aktu&#xFFFD; (*aktu&#xFFFD; (*aktu&#xFFFD; (*aktu&#xFFFD; (*aktu&#xFFFD; (*aktu&#xFFFD; (*aktu&#xFFFD; (*aktu&#xFFFD; (*aktu&#xFFFD; (*aktu&#xFFFD; (*aktu&#xFFFD; (*aktu&#xFFFD; (*aktu&#xFFFD; (*aktu&#xFFFD; (*aktu&#xFFFD; (*aktu&#xFFFD; (*aktu&#xFFFD; (*aktu&#xFFFD; (*aktu&#xFFFD; (*aktu&#xFFFD; (*aktu&#xFFFD; (*aktu&#xFFFD; (*aktu&#xFFFD; (*aktu&#xFFFD; (*aktu&#xFFFD; (*aktu&#xFFFD; (*aktu&#xFFFD; (*aktu&#xFFFD; (*aktu&#xFFFD; (*aktu&#xFFFD; (*aktu&#xFFFD; (*aktu&#xFFFD; (*aktu&#xFFFD; (*aktu&#xFFFD; (*aktu&#xFFFD; (*aktu&#xFFFD; (*aktu&#xFFFD; (*aktu&#xFFFD; (*aktu&#xFFFD; (*aktu&#xFFFD; (*aktu&#xFFFD; (*aktu&#xFFFD; (*aktu&#xFFFD; (*aktu&#xFFFD; (*aktu&#xFFFD; (*aktu&#xFFFD; (*aktu&#xFFFD; (*aktu&#xFFFD; (*aktu&#xFFFD; (*aktu&#xFFFD; (*aktu&#xFFFD; (*aktu&#xFFFD; (*aktu&#xFFFD; (*aktu&#xFFFD; (*aktu&#xFFFD; (*aktu&#xFFFD; (*aktu&#xFFFD; (*aktu&#xFFFD; (*aktu&#xFFFD; (*aktu&#xFFFD; (*aktu&#xFFFD; (*aktu&#xFFFD; (*aktu&#xFFFD; (*aktu&#xFFFD; (*aktu&#xFFFD; (*aktu&#xFFFD; (*aktu&#xFFFD; (*aktu&#xFFFD; (*aktu&#xFFFD; (*aktu&#xFFFD; (*aktu&#xFFFD; (*aktu&#xFFFD; (*aktu&#xFFFD; (*aktu&#xFFFD; (*aktu&#xFFFD; (*aktu&#xFFFD; (*aktu&#xFFFD; (*aktu&#xFFFD; (*aktu&#xFFFD; (*aktu&#xFFFD; (*aktu&#xFFFD; (*aktu&#xFFFD; (*aktu&#xFFFD; (*aktu&#xFFFD; (*aktu&#xFFFD; (*aktu&#xFFFD; (*aktu&#xFFFD; (*aktu&#xFFFD; (*aktu&#xFFFD; (*aktu&#xFFFD; (*aktu&#xFFFD; (*aktu&#xFFFD; (*aktu&#xFFFD; (*aktu&#xFFFD; (*aktu&#xFFFD; (*aktu&#xFFFD; (*aktu&#xFFFD; (*aktu&#xFFFD; (*aktu&#xFFFD; (*aktu&#xFFFD; (*aktu&#xFFFD; (*aktu&#xFFFD; (*aktu&#xFFFD; (*aktu&#xFFFD; (*aktu&#xFFFD; (*aktu&#xFFFD; (*aktu&#xFFFD; (*aktu&#xFFFD; (*aktu&#xFFFD; (*aktu&#xFFFD; (*aktu&#xFFFD; (*aktu&#xFFFD; (*aktu&#xFFFD; (*aktu&#xFFFD; (*aktu&#xFFFD; (*aktu&#xFFFD; (*aktu&#xFFFD; (*aktu&#xFFFD; (*aktu&#xFFFD; (*aktu&#xFFFD; (*aktu&#xFFFD; (*aktu&#xFFFD; (*aktu&#xFFFD; (*aktu&#xFFFD; (*aktu&#xFFFD; (*aktu&#xFFFD; (*aktu&#xFFFD; (*aktu&#xFFFD; (*aktu&#xFFFD; (*aktu&#xFFFD; (*aktu&#xFFFD; (*aktu&#xFFFD; (*aktu&#xFFFD; (*aktu&#xFFFD; (*aktu&#xFFFD; (*aktu&#xFFFD; (*aktu&#xFFFD; (*aktu&#xFFFD; (*aktu&#xFFFD; (*aktu&#xFFFD; (*aktu&#xFFFD; (*aktu&#xFFFD; (*aktu&#xFFFD; (*aktu&#xFFFD; (*aktu&#xFFFD; (*aktu&#xFFFD; (*aktu&#xFFFD; (*aktu&#xFFFD; (*aktu&#xFFFD; (*aktu&#xFFFD; (*aktu&#xFFFD; (*aktu&#xFFFD; (*aktu&#xFFFD; (*aktu&#xFFFD; (*aktu&#xFFFD; (*aktu&#xFFFD; (*aktu&#xFFFD; (*aktu&#xFFFD; (*aktu&#xFFFD; (*aktu&#xFFFD; (*aktu&#xFFFD; (*aktu&#xFFFD; (*aktu&#xFFFD; (*aktu&#xFFFD; (*aktu&#xFFFD; (*aktu&#xFFFD; (*aktu&#xFFFD; (*aktu&#xFFFD; (*aktu&#xFFFD; (*aktu&#xFFFD; (*aktu&#xFFFD; (*aktu&#xFFFD; (*aktu&#xFFFD; (*aktu&#xFFFD; (*aktu&#xFFFD; (*aktu&#xFFFD; (*aktu&#xFFFD; (*aktu&#xFFFD; (*aktu&#xFFFD; (*aktu&#xFFFD; (*aktu&#xFFFD; (*aktu&#xFFFD; (*aktu&#xFFFD; (*aktu&#xFFFD; (*aktu&#xFFFD; (*aktu&#xFFFD; (*aktu&#xFFFD; (*aktu&#xFFFD; (*aktu&#xFFFD; (*aktu&#xFFFD; (*aktu&#xFFFD; (*aktu&#xFFFD; (*aktu&#xFFFD; (*aktu&#xFFFD; (*aktu&#xFFFD; (*aktu&#xFFFD; (*aktu&#xFFFD; (*aktu&#xFFFD; (*aktu&#xFFFD; (*aktu&#xFFFD; (*aktu&#xFFFD; (*aktu&#xFFFD; (*aktu&#xFFFD; (*aktu&#xFFFD; (*aktu&#xFFFD; (*aktu&#xFFFD; (*aktu&#xFFFD; (*aktu&#xFFFD; (*aktu&#xFFFD; (*aktu&#xFFFD; (*aktu&#xFFFD; (*aktu&#xFFFD; (*aktu&#xFFFD; (*aktu&#xFFFD; (*aktu&#xFFFD; (*aktu&#xFFFD; (*aktu&#xFFFD; (*aktu&#xFFFD; (*aktu&#xFFFD; (*aktu&#xFFFD; (*aktu&#xFFFD; (*aktu&#xFFFD; (*aktu&#xFFFD; (*aktu&#xFFFD; (*aktu&#xFFFD; (*aktu&#xFFFD; (*aktu&#xFFFD; (*aktu&#xFFFD; (*aktu&#xFFFD; (*aktu&#xFFFD; (*aktu&#xFFFD; (*aktu&#xFFFD; (*aktu&#xFFFD; (*aktu&#xFFFD; (*aktu&#xFFFD; (*aktu&#xFFFD; (*aktu&#xFFFD; (*aktu&#xFFFD; (*aktu&#xFFFD; (*aktu&#xFFFD; (*aktu&#xFFFD; (*aktu&#xFFFD; (*aktu&#xFFFD; (*aktu&#xFFFD; (*aktu&#xFFFD; (*aktu&#xFFFD; (*aktu&#xFFFD; (*aktu&#xFFFD; (*aktu&#xFFFD; (*aktu&#xFFFD; (*aktu&#xFFFD; (*aktu&#xFFFD; (*aktu&#xFFFD; (*aktu&#xFFFD; (*aktu&#xFFFD; (*aktu&#xFFFD; (*aktu&#xFFFD; (*aktu&#xFFFD; (*aktu&#xFFFD; (*aktu&#xFFFD; (*aktu&#xFFFD; (*aktu&#xFFFD; (*aktu&#xFFFD; (*aktu&#xFFFD; (*aktu&#xFFFD; (*aktu&#xFFFD; (*aktu&#xFFFD; (*aktu&#xFFFD; (*aktu&#xFFFD; (*aktu&#xFFFD; (*aktu&#xFFFD; (*aktu&#xFFFD; (*aktu&#xFFFD; (*aktu&#xFFFD; (*aktu&#xFFFD; (*aktu&#xFFFD; (*aktu&#xFFFD; (*aktu&#xFFFD; (*aktu&#xFFFD; (*aktu&#xFFFD; (*aktu&#xFFFD; (*aktu&#xFFFD; (*aktu&#xFFFD; (*aktu&#xFFFD; (*aktu&#xFFFD; (*aktu&#xFFFD; (*aktu&#xFFFD; (*aktu&#xFFFD; (*aktu&#xFFFD; (*aktu&#xFFFD; (*aktu&#xFFFD; (*aktu&#xFFFD; (*aktu&#xFFFD; (*aktu&#xFFFD; (*aktu&#xFFFD; (*aktu&#xFFFD; (*aktu&#xFFFD; (*aktu&#xFFFD; (*aktu&#xFFFD; (*aktu&#xFFFD; (*aktu&#xFFFD; (*aktu&#xFFFD; (*aktu&#xFFFD; (*aktu&#xFFFD; (*aktu&#xFFFD; (*aktu&#xFFFD; (*aktu&#xFFFD; (*aktu&#xFFFD; (*aktu&#xFFFD; (*aktu&#xFFFD; (*aktu&#xFFFD; (*aktu&#xFFFD; (*aktu&#xFFFD; (*aktu&#xFFFD; (*aktu&#xFFFD; (*aktu&#xFFFD; (*aktu&#xFFFD; (*aktu&#xFFFD; (*aktu&#xFFFD; (*aktu&#xFFFD; (*aktu&#xFFFD; (*aktu&#xFFFD; (*aktu&#xFFFD; (*aktu&#xFFFD; (*aktu&#xFFFD; (*aktu&#xFFFD; (*aktu&#xFFFD; (*aktu&#xFFFD; (*aktu&#xFFFD; (*aktu&#xFFFD; (*aktu&#xFFFD; (*aktu&#xFFFD; (*aktu&#xFFFD; (*aktu&#xFFFD; (*aktu&#xFFFD; (*aktu&#xFFFD; (*aktu&#xFFFD; (*aktu&#xFFFD; (*aktu&#xFFFD; (*aktu&#xFFFD; (*aktu&#xFFFD; (*aktu&#xFFFD; (*aktu&#xFFFD; (*aktu&#xFFFD; (*aktu&#xFFFD; (*aktu&#xFFFD; (*aktu&#xFFFD; (*aktu&#xFFFD; (*aktu&#xFFFD; (*aktu&#xFFFD; (*aktu&#xFFFD; (*aktu&#xFFFD; (*aktu&#xFFFD; (*aktu&#xFFFD; (*aktu&#xFFFD; (*aktu&#xFFFD; (*aktu&#xFFFD; (*aktu&#xFFFD; (*aktu&#xFFFD; (*aktu&#xFFFD; (*aktu&#xFFFD; (*aktu&#xFFFD; (*aktu&#xFFFD; (*aktu&#xFFFD; (*aktu&#xFFFD; (*aktu&#xFFFD; (*aktu&#xFFFD; (*aktu&#xFFFD; (*aktu&#xFFFD; (*aktu&#xFFFD; (*aktu&#xFFFD; (*aktu&#xFFFD; (*aktu&#xFFFD; (*aktu&#xFFFD; (*aktu&#xFFFD; (*aktu&#xFFFD; (*aktu&#xFFFD; (*aktu&#xFFFD; (*aktu&#xFFFD; (*aktu&#xFFFD; (*aktu&#xFFFD; (*aktu&#xFFFD; (*aktu&#xFFFD; (*aktu&#xFFFD; (*aktu&#xFFFD; (*aktu&#xFFFD; (*aktu&#xFFFD; (*aktu&#xFFFD; (*aktu&#xFFFD; (*aktu&#xFFFD; (*aktu&#xFFFD; (*aktu&#xFFFD; (*aktu&#xFFFD; (*aktu&#xFFFD; (*aktu&#xFFFD; (*aktu&#xFFFD; (*aktu&#xFFFD; (*aktu&#xFFFD; (*aktu&#xFFFD; (*aktu&#xFFFD; (*aktu&#xFFFD; (*aktu&#xFFFD; (*aktu&#xFFFD; (*aktu&#xFFFD; (*aktu&#xFFFD; (*aktu&#xFFFD; (*aktu&#xFFFD; (*aktu&#xFFFD; (*aktu&#xFFFD; (*aktu&#xFFFD; (*aktu&#xFFFD; (*aktu&#xFFFD; (*aktu&#xFFFD; (*aktu&#xFFFD; (*aktu&#xFFFD; (*aktu&#xFFFD; (*aktu&#xFFFD; (*aktu&#xFFFD; (*aktu&#xFFFD; (*aktu&#xFFFD; (*aktu&#xFFFD; (*aktu&#xFFFD; (*aktu&#xFFFD; (*aktu&#xFFFD; (*aktu&#xFFFD; (*aktu&#xFFFD; (*aktu&#xFFFD; (*aktu&#xFFFD; (*aktu&#xFFFD; (*aktu&#xFFFD; (*aktu&#xFFFD; (*aktu&#xFFFD; (*aktu&#xFFFD; (*aktu&#xFFFD; (*aktu&#xFFFD; (*aktu&#xFFFD; (*aktu&#xFFFD; (*aktu&#xFFFD; (*aktu&#xFFFD; (*aktu&#xFFFD; (*aktu&#xFFFD; (*aktu&#xFFFD; (*aktu&#xFFFD; (*aktu&#xFFFD; (*aktu&#xFFFD; (*aktu&#xFFFD; (*aktu&#xFFFD; (*aktu&#xFFFD; (*aktu&#xFFFD; (*aktu&#xFFFD; (*aktu&#xFFFD; (*aktu&#xFFFD; (*aktu&#xFFFD; (*aktu&#xFFFD; (*aktu&#xFFFD; (*aktu&#xFFFD; (*aktu&#xFFFD; (*aktu&#xFFFD; (*aktu&#xFFFD; (*aktu&#xFFFD; (*aktu&#xFFFD; (*aktu&#xFFFD; (*aktu&#xFFFD; (*aktu&#xFFFD; (*aktu&#xFFFD; (*aktu&#xFFFD; (*aktu&#xFFFD; (*aktu&#xFFFD; (*aktu&#xFFFD; (*aktu&#xFFFD; (*aktu&#xFFFD; (*aktu&#xFFFD; (*aktu&#xFFFD; (*aktu&#xFFFD; (*aktu&#xFFFD; (*aktu&#xFFFD; (*aktu&#xFFFD; (*aktu&#xFFFD; (*aktu&#xFFFD; (*aktu&#xFFFD; (*aktu&#xFFFD; (*aktu&#xFFFD; (*aktu&#xFFFD; (*aktu&#xFFFD; (*aktu&#xFFFD; (*aktu&#xFFFD; (*aktu&#xFFFD; (*aktu&#xFFFD; (*aktu&#xFFFD; (*aktu&#xFFFD; (*aktu&#xFFFD; (*aktu&#xFFFD; (*aktu&#xFFFD; (*aktu&#xFFFD; (*aktu&#xFFFD; (*aktu&#xFFFD; (*aktu&#xFFFD; (*aktu&#xFFFD; (*aktu&#xFFFD; (*aktu&#xFFFD; (*aktu&#xFFFD; (*aktu&#xFFFD; (*aktu&#xFFFD; (*aktu&#xFFFD; (*aktu&#xFFFD; (*aktu&#xFFFD; (*aktu&#xFFFD; (*aktu&#xFFFD; (*aktu&#xFFFD; (*aktu&#xFFFD; (*aktu&#xFFFD; (*aktu&#xFFFD; (*aktu&#xFFFD; (*aktu&#xFFFD; (*aktu&#xFFFD; (*aktu&#xFFFD; (*aktu&#xFFFD; (*aktu&#xFFFD; (*aktu&#xFFFD; (*aktu&#xFFFD; (*aktu&#xFFFD; (*aktu&#xFFFD; (*aktu&#xFFFD; (*aktu&#xFFFD; (*aktu&#xFFFD; (*aktu&#xFFFD; (*aktu&#xFFFD; (*aktu&#xFFFD; (*aktu&#xFFFD; (*aktu&#xFFFD; (*aktu&#xFFFD; (*aktu&#xFFFD; (*aktu&#xFFFD; (*aktu&#xFFFD; (*aktu&#xFFFD; (*aktu&#xFFFD; (*aktu&#xFFFD; (*aktu&#xFFFD; (*aktu&#xFFFD; (*aktu&#xFFFD; (*aktu&#xFFFD; (*aktu&#xFFFD; (*aktu&#xFFFD; (*aktu&#xFFFD; (*aktu&#xFFFD; (*aktu&#xFFFD; (*aktu&#xFFFD; (*aktu&#xFFFD; (*aktu&#xFFFD; (*aktu&#xFFFD; (*aktu&#xFFFD; (*aktu&#xFFFD; (*aktu&#xFFFD; (*aktu&#xFFFD; (*aktu&#xFFFD; (*aktu&#xFFFD; (*aktu&#xFFFD; (*aktu&#xFFFD; (*aktu&#xFFFD; (*aktu&#xFFFD; (*aktu&#xFFFD; (*aktu&#xFFFD; (*aktu&#xFFFD; (*aktu&#xFFFD; (*aktu&#xFFFD; (*aktu&#xFFFD; (*aktu&#xFFFD; (*aktu&#xFFFD; (*aktu&#xFFFD; (*aktu&#xFFFD; (*aktu&#xFFFD; (*aktu&#xFFFD; (*aktu&#xFFFD; (*aktu&#xFFFD; (*aktu&#xFFFD; (*aktu&#xFFFD; (*aktu&#xFFFD; (*aktu&#xFFFD; (*aktu&#xFFFD; (*aktu&#xFFFD; (*aktu&#xFFFD; (*aktu&#xFFFD; (*aktu&#xFFFD; (*aktu&#xFFFD; (*aktu&#xFFFD; (*aktu&#xFFFD; (*aktu&#xFFFD; (*aktu&#xFFFD; (*aktu&#xFFFD; (*aktu&#xFFFD; (*aktu&#xFFFD; (*aktu&#xFFFD; (*aktu&#xFFFD; (*aktu&#xFFFD; (*aktu&#xFFFD; (*aktu&#xFFFD; (*aktu&#xFFFD; (*aktu&#xFFFD; (*aktu&#xFFFD; (*aktu&#xFFFD; (*aktu&#xFFFD; (*aktu&#xFFFD; (*aktu&#xFFFD; (*aktu&#xFFFD; (*aktu&#xFFFD; (*aktu&#xFFFD; (*aktu&#xFFFD; (*aktu&#xFFFD; (*aktu&#xFFFD; (*aktu&#xFFFD; (*aktu&#xFFFD; (*aktu&#xFFFD; (*aktu&#xFFFD; (*aktu&#xFFFD; (*aktu&#xFFFD; (*aktu&#xFFFD; (*aktu&#xFFFD; (*aktu&#xFFFD; (*aktu&#xFFFD; (*aktu&#xFFFD; (*aktu&#xFFFD; (*aktu&#xFFFD; (*aktu&#xFFFD; (*aktu&#xFFFD; (*aktu&#xFFFD; (*aktu&#xFFFD; (*aktu&#xFFFD; (*aktu&#xFFFD; (*aktu&#xFFFD; (*aktu&#xFFFD; (*aktu&#xFFFD; (*aktu&#xFFFD; (*aktu&#xFFFD; (*aktu&#xFFFD; (*aktu&#xFFFD; (*aktu&#xFFFD; (*aktu&#xFFFD; (*aktu&#xFFFD; (*aktu&#xFFFD; (*aktu&#xFFFD; (*aktu&#xFFFD; (*aktu&#xFFFD; (*aktu&#xFFFD; (*aktu&#xFFFD; (*aktu&#xFFFD; (*aktu&#xFFFD; (*aktu&#xFFFD; (*aktu&#xFFFD; (*aktu&#xFFFD; (*aktu&#xFFFD; (*aktu&#xFFFD; (*aktu&#xFFFD; (*aktu&#xFFFD; (*aktu&#xFFFD; (*aktu&#xFFFD; (*aktu&#xFFFD; (*aktu&#xFFFD; (*aktu&#xFFFD; (*aktu&#xFFFD; (*aktu&#xFFFD; (*aktu&#xFFFD; (*aktu&#xFFFD; (*aktu&#xFFFD; (*aktu&#xFFFD; (*aktu&#xFFFD; (*aktu&#xFFFD; (*aktu&#xFFFD; (*aktu&#xFFFD; (*aktu&#xFFFD; (*aktu&#xFFFD; (*aktu&#xFFFD; (*aktu&#xFFFD; (*aktu&#xFFFD; (*aktu&#xFFFD; (*aktu&#xFFFD; (*aktu&#xFFFD; (*aktu&#xFFFD; (*aktu&#xFFFD; (*aktu&#xFFFD; (*aktu&#xFFFD; (*aktu&#xFFFD; (*aktu&#xFFFD; (*aktu&#xFFFD; (*aktu&#xFFFD; (*aktu&#xFFFD; (*aktu&#xFFFD; (*aktu&#xFFFD; (*aktu&#xFFFD; (*aktu&#xFFFD; (*aktu&#xFFFD; (*aktu&#xFFFD; (*aktu&#xFFFD; (*aktu&#xFFFD; (*aktu&#xFFFD; (*aktu&#xFFFD; (*aktu&#xFFFD; (*aktu&#xFFFD; (*aktu&#xFFFD; (*aktu&#xFFFD; (*aktu&#xFFFD; (*aktu&#xFFFD; (*aktu&#xFFFD; (*aktu&#xFFFD; (*aktu&#xFFFD; (*aktu&#xFFFD; (*aktu&#xFFFD; (*aktu&#xFFFD; (*aktu&#xFFFD; (*aktu&#xFFFD; (*aktu&#xFFFD; (*aktu&#xFFFD; (*aktu&#xFFFD; (*aktu&#xFFFD; (*aktu&#xFFFD; (*aktu&#xFFFD; (*aktu&#xFFFD; (*aktu&#xFFFD; (*aktu&#xFFFD; (*aktu&#xFFFD; (*aktu&#xFFFD; (*aktu&#xFFFD; (*aktu&#xFFFD; (*aktu&#xFFFD; (*aktu&#xFFFD; (*aktu&#xFFFD; (*aktu&#xFFFD; (*aktu&#xFFFD; (*aktu&#xFFFD; (*aktu&#xFFFD; (*aktu&#xFFFD; (*aktu&#xFFFD; (*aktu&#xFFFD; (*aktu&#xFFFD; (*aktu&#xFFFD; (*aktu&#xFFFD; (*aktu&#xFFFD; (*aktu&#xFFFD; (*aktu&#xFFFD; (*aktu&#xFFFD; (*aktu&#xFFFD; (*aktu&#xFFFD; (*aktu&#xFFFD; (*aktu&#xFFFD; (*aktu&#xFFFD; (*aktu&#xFFFD; (*aktu&#xFFFD; (*aktu&#xFFFD; (*aktu&#xFFFD; (*aktu&#xFFFD; (*aktu&#xFFFD; (*aktu&#xFFFD; (*aktu&#xFFFD; (*aktu&#xFFFD; (*aktu&#xFFFD; (*aktu&#xFFFD; (*aktu&#xFFFD; (*aktu&#xFFFD; (*aktu&#xFFFD; (*aktu&#xFFFD; (*aktu&#xFFFD; (*aktu&#xFFFD; (*aktu&#xFFFD; (*aktu&#xFFFD; (*aktu&#xFFFD; (*aktu&#xFFFD; (*aktu&#xFFFD; (*aktu&#xFFFD; (*aktu&#xFFFD; (*aktu&#xFFFD; (*aktu&#xFFFD; (*aktu&#xFFFD; (*aktu&#xFFFD; (*aktu&#xFFFD; (*aktu&#xFFFD; (*aktu&#xFFFD; (*aktu&#xFFFD; (*aktu&#xFFFD; (*aktu&#xFFFD; (*aktu&#xFFFD; (*aktu&#xFFFD; (*aktu&#xFFFD; (*aktu&#xFFFD; (*aktu&#xFFFD; (*aktu&#xFFFD; (*aktu&#xFFFD; (*aktu&#xFFFD; (*aktu&#xFFFD; (*aktu&#xFFFD; (*aktu&#xFFFD; (*aktu&#xFFFD; (*aktu&#xFFFD; (*aktu&#xFFFD; (*aktu&#xFFFD; (*aktu&#xFFFD; (*aktu&#xFFFD; (*aktu&#xFFFD; (*aktu&#xFFFD; (*aktu&#xFFFD; (*aktu&#xFFFD; (*aktu&#xFFFD; (*aktu&#xFFFD; (*aktu&#xFFFD; (*aktu&#xFFFD; (*aktu&#xFFFD; (*aktu&#xFFFD; (*aktu&#xFFFD; (*aktu&#xFFFD; (*aktu&#xFFFD; (*aktu&#xFFFD; (*aktu&#xFFFD; (*aktu&#xFFFD; (*aktu&#xFFFD; (*aktu&#xFFFD; (*aktu&#xFFFD; (*aktu&#xFFFD; (*aktu&#xFFFD; (*aktu&#xFFFD; (*aktu&#xFFFD; (*aktu&#xFFFD; (*aktu&#xFFFD; (*aktu&#xFFFD; (*aktu&#xFFFD; (*aktu&#xFFFD; (*aktu&#xFFFD; (*aktu&#xFFFD; (*aktu&#xFFFD; (*aktu&#xFFFD; (*aktu&#xFFFD; (*aktu&#xFFFD; (*aktu&#xFFFD; (*aktu&#xFFFD; (*aktu&#xFFFD; (*aktu&#xFFFD; (*aktu&#xFFFD; (*aktu&#xFFFD; (*aktu&#xFFFD; (*aktu&#xFFFD; (*aktu&#xFFFD; (*aktu&#xFFFD; (*aktu&#xFFFD; (*aktu&#xFFFD; (*aktu&#xFFFD; (*aktu&#xFFFD; (*aktu&#xFFFD; (*aktu&#xFFFD; (*aktu&#xFFFD; (*aktu&#xFFFD; (*aktu&#xFFFD; (*aktu&#xFFFD; (*aktu&#xFFFD; (*aktu&#xFFFD; (*aktu&#xFFFD; (*aktu&#xFFFD; (*aktu&#xFFFD; (*aktu&#xFFFD; (*aktu&#xFFFD; (*aktu&#xFFFD; (*aktu&#xFFFD; (*aktu&#xFFFD; (*aktu&#xFFFD; (*aktu&#xFFFD; (*aktu&#xFFFD; (*aktu&#xFFFD; (*aktu&#xFFFD; (*aktu&#xFFFD; (*aktu&#xFFFD; (*aktu&#xFFFD; (*aktu&#xFFFD; (*aktu&#xFFFD; (*aktu&#xFFFD; (*aktu&#xFFFD; (*aktu&#xFFFD; (*aktu&#xFFFD; (*aktu&#xFFFD; (*aktu&#xFFFD; (*aktu&#xFFFD; (*aktu&#xFFFD; (*aktu&#xFFFD; (*aktu&#xFFFD; (*aktu&#xFFFD; (*aktu&#xFFFD; (*aktu&#xFFFD; (*aktu&#xFFFD; (*aktu&#xFFFD; (*aktu&#xFFFD; (*aktu&#xFFFD; (*aktu&#xFFFD; (*aktu&#xFFFD; (*aktu&#xFFFD; (*aktu&#xFFFD; (*aktu&#xFFFD; (*aktu&#xFFFD; (*aktu&#xFFFD; (*aktu&#xFFFD; (*aktu&#xFFFD; (*aktu&#xFFFD; (*aktu&#xFFFD; (*aktu&#xFFFD; (*aktu&#xFFFD; (*aktu&#xFFFD; (*aktu&#xFFFD; (*aktu&#xFFFD; (*aktu&#xFFFD; (*aktu&#xFFFD; (*aktu&#xFFFD; (*aktu&#xFFFD; (*aktu&#xFFFD; (*aktu&#xFFFD; (*aktu&#xFFFD; (*aktu&#xFFFD; (*aktu&#xFFFD; (*aktu&#xFFFD; (*aktu&#xFFFD; (*aktu&#xFFFD; (*aktu&#xFFFD; (*aktu&#xFFFD; (*aktu&#xFFFD; (*aktu&#xFFFD; (*aktu&#xFFFD; (*aktu&#xFFFD; (*aktu&#xFFFD; (*aktu&#xFFFD; (*aktu&#xFFFD; (*aktu&#xFFFD; (*aktu&#xFFFD; (*aktu&#xFFFD; (*aktu&#xFFFD; (*aktu&#xFFFD; (*aktu&#xFFFD; (*aktu&#xFFFD; (*aktu&#xFFFD; (*aktu&#xFFFD; (*aktu&#xFFFD; (*aktu&#xFFFD; (*aktu&#xFFFD; (*aktu&#xFFFD; (*aktu&#xFFFD; (*aktu&#xFFFD; (*aktu&#xFFFD; (*aktu&#xFFFD; (*aktu&#xFFFD; (*aktu&#xFFFD; (*aktu&#xFFFD; (*aktu&#xFFFD; (*aktu&#xFFFD; (*aktu&#xFFFD; (*aktu&#xFFFD; (*aktu&#xFFFD; (*aktu&#xFFFD; (*aktu&#xFFFD; (*aktu&#xFFFD; (*aktu&#xFFFD; (*aktu&#xFFFD; (*aktu&#xFFFD; (*aktu&#xFFFD; (*aktu&#xFFFD; (*aktu&#xFFFD; (*aktu&#xFFFD; (*aktu&#xFFFD; (*aktu&#xFFFD; (*aktu&#xFFFD; (*aktu&#xFFFD; (*aktu&#xFFFD; (*aktu&#xFFFD; (*aktu&#xFFFD; (*aktu&#xFFFD; (*aktu&#xFFFD; (*aktu&#xFFFD; (*aktu&#xFFFD; (*aktu&#xFFFD; (*aktu&#xFFFD; (*aktu&#xFFFD; (*aktu&#xFFFD; (*aktu&#xFFFD; (*aktu&#xFFFD; (*aktu&#xFFFD; (*aktu&#xFFFD; (*aktu&#xFFFD; (*aktu&#xFFFD; (*aktu&#xFFFD; (*aktu&#xFFFD; (*aktu&#xFFFD; (*aktu&#xFFFD; (*aktu&#xFFFD; (*aktu&#xFFFD; (*aktu&#xFFFD; (*aktu&#xFFFD; (*aktu&#xFFFD; (*aktu&#xFFFD; (*aktu&#xFFFD; (*aktu&#xFFFD; (*aktu&#xFFFD; (*aktu&#xFFFD; (*aktu&#xFFFD; (*aktu&#xFFFD; (*aktu&#xFFFD; (*aktu&#xFFFD; (*aktu&#xFFFD; (*aktu&#xFFFD; (*aktu&#xFFFD; (*aktu&#xFFFD; (*aktu&#xFFFD; (*aktu&#xFFFD; (*aktu&#xFFFD; (*aktu&#xFFFD; (*aktu&#xFFFD; (*aktu&#xFFFD; (*aktu&#xFFFD; (*aktu&#xFFFD; (*aktu&#xFFFD; (*aktu&#xFFFD; (*aktu&#xFFFD; (*aktu&#xFFFD; (*aktu&#xFFFD; (*aktu&#xFFFD; (*aktu&#xFFFD; (*aktu&#xFFFD; (*aktu&#xFFFD; (*aktu&#xFFFD; (*aktu&#xFFFD; (*aktu&#xFFFD; (*aktu&#xFFFD; (*aktu&#xFFFD; (*aktu&#xFFFD; (*aktu&#xFFFD; (*aktu&#xFFFD; (*aktu&#xFFFD; (*aktu&#xFFFD; (*aktu&#xFFFD; (*aktu&#xFFFD; (*aktu&#xFFFD; (*aktu&#xFFFD; (*aktu&#xFFFD; (*aktu&#xFFFD; (*aktu&#xFFFD; (*aktu&#xFFFD; (*aktu&#xFFFD; (*aktu&#xFFFD; (*aktu&#xFFFD; (*aktu&#xFFFD; (*aktu&#xFFFD; (*aktu&#xFFFD; (*aktu&#xFFFD; (*aktu&#xFFFD; (*aktu&#xFFFD; (*aktu&#xFFFD; (*aktu&#xFFFD; (*aktu&#xFFFD; (*aktu&#xFFFD; (*aktu&#xFFFD; (*aktu&#xFFFD; (*aktu&#xFFFD; (*aktu&#xFFFD; (*aktu&#xFFFD; (*aktu&#xFFFD; (*aktu&#xFFFD; (*aktu&#xFFFD; (*aktu&#xFFFD; (*aktu&#xFFFD; (*aktu&#xFFFD; (*aktu&#xFFFD; (*aktu&#xFFFD; (*aktu&#xFFFD; (*aktu&#xFFFD; (*aktu&#xFFFD; (*aktu&#xFFFD; (*aktu&#xFFFD; (*aktu&#xFFFD; (*aktu&#xFFFD; (*aktu&#xFFFD; (*aktu&#xFFFD; (*aktu&#xFFFD; (*aktu&#xFFFD; (*aktu&#xFFFD; (*aktu&#xFFFD; (*aktu&#xFFFD; (*aktu&#xFFFD; (*aktu&#xFFFD; (*aktu&#xFFFD; (*aktu&#xFFFD; (*aktu&#xFFFD; (*aktu&#xFFFD; (*aktu&#xFFFD; (*aktu&#xFFFD; (*aktu&#xFFFD; (*aktu&#xFFFD; (*aktu&#xFFFD; (*aktu&#xFFFD; (*aktu&#xFFFD; (*aktu&#xFFFD; (*aktu&#xFFFD; (*aktu&#xFFFD; (*aktu&#xFFFD; (*aktu&#xFFFD; (*aktu&#xFFFD; (*aktu&#xFFFD; (*aktu&#xFFFD; (*aktu&#xFFFD; (*aktu&#xFFFD; (*aktu&#xFFFD; (*aktu&#xFFFD; (*aktu&#xFFFD; (*aktu&#xFFFD; (*aktu&#xFFFD; (*aktu&#xFFFD; (*aktu&#xFFFD; (*aktu&#xFFFD; (*aktu&#xFFFD; (*aktu&#xFFFD; (*aktu&#xFFFD; (*aktu&#xFFFD; (*aktu&#xFFFD; (*aktu&#xFFFD; (*aktu&#xFFFD; (*aktu&#xFFFD; (*aktu&#xFFFD; (*aktu&#xFFFD; (*aktu&#xFFFD; (*aktu&#xFFFD; (*aktu&#xFFFD; (*aktu&#xFFFD; (*aktu&#xFFFD; (*aktu&#xFFFD; (*aktu&#xFFFD; (*aktu&#xFFFD; (*aktu&#xFFFD; (*aktu&#xFFFD; (*aktu&#xFFFD; (*aktu&#xFFFD; (*aktu&#xFFFD; (*aktu&#xFFFD; (*aktu&#xFFFD; (*aktu&#xFFFD; (*aktu&#xFFFD; (*aktu&#xFFFD; (*aktu&#xFFFD; (*aktu&#xFFFD; (*aktu&#xFFFD; (*aktu&#xFFFD; (*aktu&#xFFFD; (*aktu&#xFFFD; (*aktu&#xFFFD; (*aktu&#xFFFD; (*aktu&#xFFFD; (*aktu&#xFFFD; (*aktu&#xFFFD; (*aktu&#xFFFD; (*aktu&#xFFFD; (*aktu&#xFFFD; (*aktu&#xFFFD; (*aktu&#xFFFD; (*aktu&#xFFFD; (*aktu&#xFFFD; (*aktu&#xFFFD; (*aktu&#xFFFD; (*aktu&#xFFFD; (*aktu&#xFFFD; (*aktu&#xFFFD; (*aktu&#xFFFD; (*aktu&#xFFFD; (*aktu&#xFFFD; (*aktu&#xFFFD; (*aktu&#xFFFD; (*aktu&#xFFFD; (*aktu&#xFFFD; (*aktu&#xFFFD; (*aktu&#xFFFD; (*aktu&#xFFFD; (*aktu&#xFFFD; (*aktu&#xFFFD; (*aktu&#xFFFD; (*aktu&#xFFFD; (*aktu&#xFFFD; (*aktu&#xFFFD; (*aktu&#xFFFD; (*aktu&#xFFFD; (*aktu&#xFFFD; (*aktu&#xFFFD; (*aktu&#xFFFD; (*aktu&#xFFFD; (*aktu&#xFFFD; (*aktu&#xFFFD; (*aktu&#xFFFD; (*aktu&#xFFFD; (*aktu&#xFFFD; (*aktu&#xFFFD; (*aktu&#xFFFD; (*aktu&#xFFFD; (*aktu&#xFFFD; (*aktu&#xFFFD; (*aktu&#xFFFD; (*aktu&#xFFFD; (*aktu&#xFFFD; (*aktu&#xFFFD; (*aktu&#xFFFD; (*aktu&#xFFFD; (*aktu&#xFFFD; (*aktu&#xFFFD; (*aktu&#xFFFD; (*aktu&#xFFFD; (*aktu&#xFFFD; (*aktu&#xFFFD; (*aktu&#xFFFD; (*aktu&#xFFFD; (*aktu&#xFFFD; (*aktu&#xFFFD; (*aktu&#xFFFD; (*aktu&#xFFFD; (*aktu&#xFFFD; (*aktu&#xFFFD; (*aktu&#xFFFD; (*aktu&#xFFFD; (*aktu&#xFFFD; (*aktu&#xFFFD; (*aktu&#xFFFD; (*aktu&#xFFFD; (*aktu&#xFFFD; (*aktu&#xFFFD; (*aktu&#xFFFD; (*aktu&#xFFFD; (*aktu&#xFFFD; (*aktu&#xFFFD; (*aktu&#xFFFD; (*aktu&#xFFFD; (*aktu&#xFFFD; (*aktu&#xFFFD; (*aktu&#xFFFD; (*aktu&#xFFFD; (*aktu&#xFFFD; (*aktu&#xFFFD; (*aktu&#xFFFD; (*aktu&#xFFFD; (*aktu&#xFFFD; (*aktu&#xFFFD; (*aktu&#xFFFD; (*aktu&#xFFFD; (*aktu&#xFFFD; (*aktu&#xFFFD; (*aktu&#xFFFD; (*aktu&#xFFFD; (*aktu&#xFFFD; (*aktu&#xFFFD; (*aktu&#xFFFD; (*aktu&#xFFFD; (*aktu&#xFFFD; (*aktu&#xFFFD; (*aktu&#xFFFD; (*aktu&#xFFFD; (*aktu&#xFFFD; (*aktu&#xFFFD; (*aktu&#xFFFD; (*aktu&#xFFFD; (*aktu&#xFFFD; (*aktu&#xFFFD; (*aktu&#xFFFD; (*aktu&#xFFFD; (*aktu&#xFFFD; (*aktu&#xFFFD; (*aktu&#xFFFD; (*aktu&#xFFFD; (*aktu&#xFFFD; (*aktu&#xFFFD; (*aktu&#xFFFD; (*aktu&#xFFFD; (*aktu&#xFFFD; (*aktu&#xFFFD; (*aktu&#xFFFD; (*aktu&#xFFFD; (*aktu&#xFFFD; (*aktu&#xFFFD; (*aktu&#xFFFD; (*aktu&#xFFFD; (*aktu&#xFFFD; (*aktu&#xFFFD; (*aktu&#xFFFD; (*aktu&#xFFFD; (*aktu&#xFFFD; (*aktu&#xFFFD; (*aktu&#xFFFD; (*aktu&#xFFFD; (*aktu&#xFFFD; (*aktu&#xFFFD; (*aktu&#xFFFD; (*aktu&#xFFFD; (*aktu&#xFFFD; (*aktu&#xFFFD; (*aktu&#xFFFD; (*aktu&#xFFFD; (*aktu&#xFFFD; (*aktu&#xFFFD; (*aktu&#xFFFD; (*aktu&#xFFFD; (*aktu&#xFFFD; (*aktu&#xFFFD; (*aktu&#xFFFD; (*aktu&#xFFFD; (*aktu&#xFFFD; (*aktu&#xFFFD; (*aktu&#xFFFD; (*aktu&#xFFFD; (*aktu&#xFFFD; (*aktu&#xFFFD; (*aktu&#xFFFD; (*aktu&#xFFFD; (*aktu&#xFFFD; (*aktu&#xFFFD; (*aktu&#xFFFD; (*aktu&#xFFFD; (*aktu&#xFFFD; (*aktu&#xFFFD; (*aktu&#xFFFD; (*aktu&#xFFFD; (*aktu&#xFFFD; (*aktu&#xFFFD; (*aktu&#xFFFD; (*aktu&#xFFFD; (*aktu&#xFFFD; (*aktu&#xFFFD; (*aktu&#xFFFD; (*aktu&#xFFFD; (*aktu&#xFFFD; (*aktu&#xFFFD; (*aktu&#xFFFD; (*aktu&#xFFFD; (*aktu&#xFFFD; (*aktu&#xFFFD; (*aktu&#xFFFD; (*aktu&#xFFFD; (*aktu&#xFFFD; (*aktu&#xFFFD; (*aktu&#xFFFD; (*aktu&#xFFFD; (*aktu&#xFFFD; (*aktu&#xFFFD; (*aktu&#xFFFD; (*aktu&#xFFFD; (*aktu&#xFFFD; (*aktu&#xFFFD; (*aktu&#xFFFD; (*aktu&#xFFFD; (*aktu&#xFFFD; (*aktu&#xFFFD; (*aktu&#xFFFD; (*aktu&#xFFFD; (*aktu&#xFFFD; (*aktu&#xFFFD; (*aktu&#xFFFD; (*aktu&#xFFFD; (*aktu&#xFFFD; (*aktu&#xFFFD; (*aktu&#xFFFD; (*aktu&#xFFFD; (*aktu&#xFFFD; (*aktu&#xFFFD; (*aktu&#xFFFD; (*aktu&#xFFFD; (*aktu&#xFFFD; (*aktu&#xFFFD; (*aktu&#xFFFD; (*aktu&#xFFFD; (*aktu&#xFFFD; (*aktu&#xFFFD; (*aktu&#xFFFD; (*aktu&#xFFFD; (*aktu&#xFFFD; (*aktu&#xFFFD; (*aktu&#xFFFD; (*aktu&#xFFFD; (*aktu&#xFFFD; (*aktu&#xFFFD; (*aktu&#xFFFD; (*aktu&#xFFFD; (*aktu&#xFFFD; (*aktu&#xFFFD; (*aktu&#xFFFD; (*aktu&#xFFFD; (*aktu&#xFFFD; (*aktu&#xFFFD; (*aktu&#xFFFD; (*aktu&#xFFFD; (*aktu&#xFFFD; (*aktu&#xFFFD; (*aktu&#xFFFD; (*aktu&#xFFFD; (*aktu&#xFFFD; (*aktu&#xFFFD; (*aktu&#xFFFD; (*aktu&#xFFFD; (*aktu&#xFFFD; (*aktu&#xFFFD; (*aktu&#xFFFD; (*aktu&#xFFFD; (*aktu&#xFFFD; (*aktu&#xFFFD; (*aktu&#xFFFD; (*aktu&#xFFFD; (*aktu&#xFFFD; (*aktu&#xFFFD; (*aktu&#xFFFD; (*aktu&#xFFFD; (*aktu&#xFFFD; (*aktu&#xFFFD; (*aktu&#xFFFD; (*aktu&#xFFFD; (*aktu&#xFFFD; (*aktu&#xFFFD; (*aktu&#xFFFD; (*aktu&#xFFFD; (*aktu&#xFFFD; (*aktu&#xFFFD; (*aktu&#xFFFD; (*aktu&#xFFFD; (*aktu&#xFFFD; (*aktu&#xFFFD; (*aktu&#xFFFD; (*aktu&#xFFFD; (*aktu&#xFFFD; (*aktu&#xFFFD; (*aktu&#xFFFD; (*aktu&#xFFFD; (*aktu&#xFFFD; (*aktu&#xFFFD; (*aktu&#xFFFD; (*aktu&#xFFFD; (*aktu&#xFFFD; (*aktu&#xFFFD; (*aktu&#xFFFD; (*aktu&#xFFFD; (*aktu&#xFFFD; (*aktu&#xFFFD; (*aktu&#xFFFD; (*aktu&#xFFFD; (*aktu&#xFFFD; (*aktu&#xFFFD; (*aktu&#xFFFD; (*aktu&#xFFFD; (*aktu&#xFFFD; (*aktu&#xFFFD; (*aktu&#xFFFD; (*aktu&#xFFFD; (*aktu&#xFFFD; (*aktu&#xFFFD; (*aktu&#xFFFD; (*aktu&#xFFFD; (*aktu&#xFFFD; (*aktu&#xFFFD; (*aktu&#xFFFD; (*aktu&#xFFFD; (*aktu&#xFFFD; (*aktu&#xFFFD; (*aktu&#xFFFD; (*aktu&#xFFFD; (*aktu&#xFFFD; (*aktu&#xFFFD; (*aktu&#xFFFD; (*aktu&#xFFFD; (*aktu&#xFFFD; (*aktu&#xFFFD; (*aktu&#xFFFD; (*aktu&#xFFFD; (*aktu&#xFFFD; (*aktu&#xFFFD; (*aktu&#xFFFD; (*aktu&#xFFFD; (*aktu&#xFFFD; (*aktu&#xFFFD; (*aktu&#xFFFD; (*aktu&#xFFFD; (*aktu&#xFFFD; (*aktu&#xFFFD; (*aktu&#xFFFD; (*aktu&#xFFFD; (*aktu&#xFFFD; (*aktu&#xFFFD; (*aktu&#xFFFD; (*aktu&#xFFFD; (*aktu&#xFFFD; (*aktu&#xFFFD; (*aktu&#xFFFD; (*aktu&#xFFFD; (*aktu&#xFFFD; (*aktu&#xFFFD; (*aktu&#xFFFD; (*aktu&#xFFFD; (*aktu&#xFFFD; (*aktu&#xFFFD; (*aktu&#xFFFD; (*aktu&#xFFFD; (*aktu&#xFFFD; (*aktu&#xFFFD; (*aktu&#xFFFD; (*aktu&#xFFFD; (*aktu&#xFFFD; (*aktu&#xFFFD; (*aktu&#xFFFD; (*aktu&#xFFFD; (*aktu&#xFFFD; (*aktu&#xFFFD; (*aktu&#xFFFD; (*aktu&#xFFFD; (*aktu&#xFFFD; (*aktu&#xFFFD; (*aktu&#xFFFD; (*aktu&#xFFFD; (*aktu&#xFFFD; (*aktu&#xFFFD; (*aktu&#xFFFD; (*aktu&#xFFFD; (*aktu&#xFFFD; (*aktu&#xFFFD; (*aktu&#xFFFD; (*aktu&#xFFFD; (*aktu&#xFFFD; (*aktu&#xFFFD; (*aktu&#xFFFD; (*aktu&#xFFFD; (*aktu&#xFFFD; (*aktu&#xFFFD; (*aktu&#xFFFD; (*aktu&#xFFFD; (*aktu&#xFFFD; (*aktu&#xFFFD; (*aktu&#xFFFD; (*aktu&#xFFFD; (*aktu&#xFFFD; (*aktu&#xFFFD; (*aktu&#xFFFD; (*aktu&#xFFFD; (*aktu&#xFFFD; (*aktu&#xFFFD; (*aktu&#xFFFD; (*aktu&#xFFFD; (*aktu&#xFFFD; (*aktu&#xFFFD; (*aktu&#xFFFD; (*aktu&#xFFFD; (*aktu&#xFFFD; (*aktu&#xFFFD; (*aktu&#xFFFD; (*aktu&#xFFFD; (*aktu&#xFFFD; (*aktu&#xFFFD; (*aktu&#xFFFD; (*aktu&#xFFFD; (*aktu&#xFFFD; (*aktu&#xFFFD; (*aktu&#xFFFD; (*aktu&#xFFFD; (*aktu&#xFFFD; (*aktu&#xFFFD; (*aktu&#xFFFD; (*aktu&#xFFFD; (*aktu&#xFFFD; (*aktu&#xFFFD; (*aktu&#xFFFD; (*aktu&#xFFFD; (*aktu&#xFFFD; (*aktu&#xFFFD; (*aktu&#xFFFD; (*aktu&#xFFFD; (*aktu&#xFFFD; (*aktu&#xFFFD; (*aktu&#xFFFD; (*aktu&#xFFFD; (*aktu&#xFFFD; (*aktu&#xFFFD; (*aktu&#xFFFD; (*aktu&#xFFFD; (*aktu&#xFFFD; (*aktu&#xFFFD; (*aktu&#xFFFD; (*aktu&#xFFFD; (*aktu&#xFFFD; (*aktu&#xFFFD; (*aktu&#xFFFD; (*aktu&#xFFFD; (*aktu&#xFFFD; (*aktu&#xFFFD; (*aktu&#xFFFD; (*aktu&#xFFFD; (*aktu&#xFFFD; (*aktu&#xFFFD; (*aktu&#xFFFD; (*aktu&#xFFFD; (*aktu&#xFFFD; (*aktu&#xFFFD; (*aktu&#xFFFD; (*aktu&#xFFFD; (*aktu&#xFFFD; (*aktu&#xFFFD; (*aktu&#xFFFD; (*aktu&#xFFFD; (*aktu&#xFFFD; (*aktu&#xFFFD; (*aktu&#xFFFD; (*aktu&#xFFFD; (*aktu&#xFFFD; (*aktu&#xFFFD; (*aktu&#xFFFD; (*aktu&#xFFFD; (*aktu&#xFFFD; (*aktu&#xFFFD; (*aktu&#xFFFD; (*aktu&#xFFFD; (*aktu&#xFFFD; (*aktu&#xFFFD; (*aktu&#xFFFD; (*aktu&#xFFFD; (*aktu&#xFFFD; (*aktu&#xFFFD; (*aktu&#xFFFD; (*aktu&#xFFFD; (*aktu&#xFFFD; (*aktu&#xFFFD; (*aktu&#xFFFD; (*aktu&#xFFFD; (*aktu&#xFFFD; (*aktu&#xFFFD; (*aktu&#xFFFD; (*aktu&#xFFFD; (*aktu&#xFFFD; (*aktu&#xFFFD; (*aktu&#xFFFD; (*aktu&#xFFFD; (*aktu&#xFFFD; (*aktu&#xFFFD; (*aktu&#xFFFD; (*aktu&#xFFFD; (*aktu&#xFFFD; (*aktu&#xFFFD; (*aktu&#xFFFD; (*aktu&#xFFFD; (*aktu&#xFFFD; (*aktu&#xFFFD; (*aktu&#xFFFD; (*aktu&#xFFFD; (*aktu&#xFFFD; (*aktu&#xFFFD; (*aktu&#xFFFD; (*aktu&#xFFFD; (*aktu&#xFFFD; (*aktu&#xFFFD; (*aktu&#xFFFD; (*aktu&#xFFFD; (*aktu&#xFFFD; (*aktu&#xFFFD; (*aktu&#xFFFD; (*aktu&#xFFFD; (*aktu&#xFFFD; (*aktu&#xFFFD; (*aktu&#xFFFD; (*aktu&#xFFFD; (*aktu&#xFFFD; (*aktu&#xFFFD; (*aktu&#xFFFD; (*aktu&#xFFFD; (*aktu&#xFFFD; (*aktu&#xFFFD; (*aktu&#xFFFD; (*aktu&#xFFFD; (*aktu&#xFFFD; (*aktu&#xFFFD; (*aktu&#xFFFD; (*aktu&#xFFFD; (*aktu&#xFFFD; (*aktu&#xFFFD; (*aktu&#xFFFD; (*aktu&#xFFFD; (*aktu&#xFFFD; (*aktu&#xFFFD; (*aktu&#xFFFD; (*aktu&#xFFFD; (*aktu&#xFFFD; (*aktu&#xFFFD; (*aktu&#xFFFD; (*aktu&#xFFFD; (*aktu&#xFFFD; (*aktu&#xFFFD; (*aktu&#xFFFD; (*aktu&#xFFFD; (*aktu&#xFFFD; (*aktu&#xFFFD; (*aktu&#xFFFD; (*aktu&#xFFFD; (*aktu&#xFFFD; (*aktu&#xFFFD; (*aktu&#xFFFD; (*aktu&#xFFFD; (*aktu&#xFFFD; (*aktu&#xFFFD; (*aktu&#xFFFD; (*aktu&#xFFFD; (*aktu&#xFFFD; (*aktu&#xFFFD; (*aktu&#xFFFD; (*aktu&#xFFFD; (*aktu&#xFFFD; (*aktu&#xFFFD; (*aktu&#xFFFD; (*aktu&#xFFFD; (*aktu&#xFFFD; (*aktu&#xFFFD; (*aktu&#xFFFD; (*aktu&#xFFFD; (*aktu&#xFFFD; (*aktu&#xFFFD; (*aktu&#xFFFD; (*aktu&#xFFFD; (*aktu&#xFFFD; (*aktu&#xFFFD; (*aktu&#xFFFD; (*aktu&#xFFFD; (*aktu&#xFFFD; (*aktu&#xFFFD; (*aktu&#xFFFD; (*aktu&#xFFFD; (*aktu&#xFFFD; (*aktu&#xFFFD; (*aktu&#xFFFD; (*aktu&#xFFFD; (*aktu&#xFFFD; (*aktu&#xFFFD; (*aktu&#xFFFD; (*aktu&#xFFFD; (*aktu&#xFFFD; (*aktu&#xFFFD; (*aktu&#xFFFD; (*aktu&#xFFFD; (*aktu&#xFFFD; (*aktu&#xFFFD; (*aktu&#xFFFD; (*aktu&#xFFFD; (*aktu&#xFFFD; (*aktu&#xFFFD; (*aktu&#xFFFD; (*aktu&#xFFFD; (*aktu&#xFFFD; (*aktu&#xFFFD; (*aktu&#xFFFD; (*aktu&#xFFFD; (*aktu&#xFFFD; (*aktu&#xFFFD; (*aktu&#xFFFD; (*aktu&#xFFFD; (*aktu&#xFFFD; (*aktu&#xFFFD; (*aktu&#xFFFD; (*aktu&#xFFFD; (*aktu&#xFFFD; (*aktu&#xFFFD; (*aktu&#xFFFD; (*aktu&#xFFFD; (*aktu&#xFFFD; (*aktu&#xFFFD; (*aktu&#xFFFD; (*aktu&#xFFFD; (*aktu&#xFFFD; (*aktu&#xFFFD; (*aktu&#xFFFD; (*aktu&#xFFFD; (*aktu&#xFFFD; (*aktu&#xFFFD; (*aktu&#xFFFD; (*aktu&#xFFFD; (*aktu&#xFFFD; (*aktu&#xFFFD; (*aktu&#xFFFD; (*aktu&#xFFFD; (*aktu&#xFFFD; (*aktu&#xFFFD; (*aktu&#xFFFD; (*aktu&#xFFFD; (*aktu&#xFFFD; (*aktu&#xFFFD; (*aktu&#xFFFD; (*aktu&#xFFFD; (*aktu&#xFFFD; (*aktu&#xFFFD; (*aktu&#xFFFD; (*aktu&#xFFFD; (*aktu&#xFFFD; (*aktu&#xFFFD; (*aktu&#xFFFD; (*aktu&#xFFFD; (*aktu&#xFFFD; (*aktu&#xFFFD; (*aktu&#xFFFD; (*aktu&#xFFFD; (*aktu&#xFFFD; (*aktu&#xFFFD; (*aktu&#xFFFD; (*aktu&#xFFFD; (*aktu&#xFFFD; (*aktu&#xFFFD; (*aktu&#xFFFD; (*aktu&#xFFFD; (*aktu&#xFFFD; (*aktu&#xFFFD; (*aktu&#xFFFD; (*aktu&#xFFFD; (*aktu&#xFFFD; (*aktu&#xFFFD; (*aktu&#xFFFD; (*aktu&#xFFFD; (*aktu&#xFFFD; (*aktu&#xFFFD; (*aktu&#xFFFD; (*aktu&#xFFFD; (*aktu&#xFFFD; (*aktu&#xFFFD; (*aktu&#xFFFD; (*aktu&#xFFFD; (*aktu&#xFFFD; (*aktu&#xFFFD; (*aktu&#xFFFD; (*aktu&#xFFFD; (*aktu&#xFFFD; (*aktu&#xFFFD; (*aktu&#xFFFD; (*aktu&#xFFFD; (*aktu&#xFFFD; (*aktu&#xFFFD; (*aktu&#xFFFD; (*aktu&#xFFFD; (*aktu&#xFFFD; (*aktu&#xFFFD; (*aktu&#xFFFD; (*aktu&#xFFFD; (*aktu&#xFFFD; (*aktu&#xFFFD; (*aktu&#xFFFD; (*aktu&#xFFFD; (*aktu&#xFFFD; (*aktu&#xFFFD; (*aktu&#xFFFD; (*aktu&#xFFFD; (*aktu&#xFFFD; (*aktu&#xFFFD; (*aktu&#xFFFD; (*aktu&#xFFFD; (*aktu&#xFFFD; (*aktu&#xFFFD; (*aktu&#xFFFD; (*aktu&#xFFFD; (*aktu&#xFFFD; (*aktu&#xFFFD; (*aktu&#xFFFD; (*aktu&#xFFFD; (*aktu&#xFFFD; (*aktu&#xFFFD; (*aktu&#xFFFD; (*aktu&#xFFFD; (*aktu&#xFFFD; (*aktu&#xFFFD; (*aktu&#xFFFD; (*aktu&#xFFFD; (*aktu&#xFFFD; (*aktu&#xFFFD; (*aktu&#xFFFD; (*aktu&#xFFFD; (*aktu&#xFFFD; (*aktu&#xFFFD; (*aktu&#xFFFD; (*aktu&#xFFFD; (*aktu&#xFFFD; (*aktu&#xFFFD; (*aktu&#xFFFD; (*aktu&#xFFFD; (*aktu&#xFFFD; (*aktu&#xFFFD; (*aktu&#xFFFD; (*aktu&#xFFFD; (*aktu&#xFFFD; (*aktu&#xFFFD; (*aktu&#xFFFD; (*aktu&#xFFFD; (*aktu&#xFFFD; (*aktu&#xFFFD; (*aktu&#xFFFD; (*aktu&#xFFFD; (*aktu&#xFFFD; (*aktu&#xFFFD; (*aktu&#xFFFD; (*aktu&#xFFFD; (*aktu&#xFFFD; (*aktu&#xFFFD; (*aktu&#xFFFD; (*aktu&#xFFFD; (*aktu&#xFFFD; (*aktu&#xFFFD; (*aktu&#xFFFD; (*aktu&#xFFFD; (*aktu&#xFFFD; (*aktu&#xFFFD; (*aktu&#xFFFD; (*aktu&#xFFFD; (*aktu&#xFFFD; (*aktu&#xFFFD; (*aktu&#xFFFD; (*aktu&#xFFFD; (*aktu&#xFFFD; (*aktu&#xFFFD; (*aktu&#xFFFD; (*aktu&#xFFFD; (*aktu&#xFFFD; (*aktu&#xFFFD; (*aktu&#xFFFD; (*aktu&#xFFFD; (*aktu&#xFFFD; (*aktu&#xFFFD; (*aktu&#xFFFD; (*aktu&#xFFFD; (*aktu&#xFFFD; (*aktu&#xFFFD; (*aktu&#xFFFD; (*aktu&#xFFFD; (*aktu&#xFFFD; (*aktu&#xFFFD; (*aktu&#xFFFD; (*aktu&#xFFFD; (*aktu&#xFFFD; (*aktu&#xFFFD; (*aktu&#xFFFD; (*aktu&#xFFFD; (*aktu&#xFFFD; (*aktu&#xFFFD; (*aktu&#xFFFD; (*aktu&#xFFFD; (*aktu&#xFFFD; (*aktu&#xFFFD; (*aktu&#xFFFD; (*aktu&#xFFFD; (*aktu&#xFFFD; (*aktu&#xFFFD; (*aktu&#xFFFD; (*aktu&#xFFFD; (*aktu&#xFFFD; (*aktu&#xFFFD; (*aktu&#xFFFD; (*aktu&#xFFFD; (*aktu&#xFFFD; (*aktu&#xFFFD; (*aktu&#xFFFD; (*aktu&#xFFFD; (*aktu&#xFFFD; (*aktu&#xFFFD; (*aktu&#xFFFD; (*aktu&#xFFFD; (*aktu&#xFFFD; (*aktu&#xFFFD; (*aktu&#xFFFD; (*aktu&#xFFFD; (*aktu&#xFFFD; (*aktu&#xFFFD; (*aktu&#xFFFD; (*aktu&#xFFFD; (*aktu&#xFFFD; (*aktu&#xFFFD; (*aktu&#xFFFD; (*aktu&#xFFFD; (*aktu&#xFFFD; (*aktu&#xFFFD; (*aktu&#xFFFD; (*aktu&#xFFFD; (*aktu&#xFFFD; (*aktu&#xFFFD; (*aktu&#xFFFD; (*aktu&#xFFFD; (*aktu&#xFFFD; (*aktu&#xFFFD; (*aktu&#xFFFD; (*aktu&#xFFFD; (*aktu&#xFFFD; (*aktu&#xFFFD; (*aktu&#xFFFD; (*aktu&#xFFFD; (*aktu&#xFFFD; (*aktu&#xFFFD; (*aktu&#xFFFD; (*aktu&#xFFFD; (*aktu&#xFFFD; (*aktu&#xFFFD; (*aktu&#xFFFD; (*aktu&#xFFFD; (*aktu&#xFFFD; (*aktu&#xFFFD; (*aktu&#xFFFD; (*aktu&#xFFFD; (*aktu&#xFFFD; (*aktu&#xFFFD; (*aktu&#xFFFD; (*aktu&#xFFFD; (*aktu&#xFFFD; (*aktu&#xFFFD; (*aktu&#xFFFD; (*aktu&#xFFFD; (*aktu&#xFFFD; (*aktu&#xFFFD; (*aktu&#xFFFD; (*aktu&#xFFFD; (*aktu&#xFFFD; (*aktu&#xFFFD; (*aktu&#xFFFD; (*aktu&#xFFFD; (*aktu&#xFFFD; (*aktu&#xFFFD; (*aktu&#xFFFD; (*aktu&#xFFFD; (*aktu&#xFFFD; (*aktu&#xFFFD; (*aktu&#xFFFD; (*aktu&#xFFFD; (*aktu&#xFFFD; (*aktu&#xFFFD; (*aktu&#xFFFD; (*aktu&#xFFFD; (*aktu&#xFFFD; (*aktu&#xFFFD; (*aktu&#xFFFD; (*aktu&#xFFFD; (*aktu&#xFFFD; (*aktu&#xFFFD; (*aktu&#xFFFD; (*aktu&#xFFFD; (*aktu&#xFFFD; (*aktu&#xFFFD; (*aktu&#xFFFD; (*aktu&#xFFFD; (*aktu&#xFFFD; (*aktu&#xFFFD; (*aktu&#xFFFD; (*aktu&#xFFFD; (*aktu&#xFFFD; (*aktu&#xFFFD; (*aktu&#xFFFD; (*aktu&#xFFFD; (*aktu&#xFFFD; (*aktu&#xFFFD; (*aktu&#xFFFD; (*aktu&#xFFFD; (*aktu&#xFFFD; (*aktu&#xFFFD; (*aktu&#xFFFD; (*aktu&#xFFFD; (*aktu&#xFFFD; (*aktu&#xFFFD; (*aktu&#xFFFD; (*aktu&#xFFFD; (*aktu&#xFFFD; (*aktu&#xFFFD; (*aktu&#xFFFD; (*aktu&#xFFFD; (*aktu&#xFFFD; (*aktu&#xFFFD; (*aktu&#xFFFD; (*aktu&#xFFFD; (*aktu&#xFFFD; (*aktu&#xFFFD; (*aktu&#xFFFD; (*aktu&#xFFFD; (*aktu&#xFFFD; (*aktu&#xFFFD; (*aktu&#xFFFD; (*aktu&#xFFFD; (*aktu&#xFFFD; (*aktu&#xFFFD; (*aktu&#xFFFD; (*aktu&#xFFFD; (*aktu&#xFFFD; (*aktu&#xFFFD; (*aktu&#xFFFD; (*aktu&#xFFFD; (*aktu&#xFFFD; (*aktu&#xFFFD; (*aktu&#xFFFD; (*aktu&#xFFFD; (*aktu&#xFFFD; (*aktu&#xFFFD; (*aktu&#xFFFD; (*aktu&#xFFFD; (*aktu&#xFFFD; (*aktu&#xFFFD; (*aktu&#xFFFD; (*aktu&#xFFFD; (*aktu&#xFFFD; (*aktu&#xFFFD; (*aktu&#xFFFD; (*aktu&#xFFFD; (*aktu&#xFFFD; (*aktu&#xFFFD; (*aktu&#xFFFD; (*aktu&#xFFFD; (*aktu&#xFFFD; (*aktu&#xFFFD; (*aktu&#xFFFD; (*aktu&#xFFFD; (*aktu&#xFFFD; (*aktu&#xFFFD; (*aktu&#xFFFD; (*aktu&#xFFFD; (*aktu&#xFFFD; (*aktu&#xFFFD; (*aktu&#xFFFD; (*aktu&#xFFFD; (*aktu&#xFFFD; (*aktu&#xFFFD; (*aktu&#xFFFD; (*aktu&#xFFFD; (*aktu&#xFFFD; (*aktu&#xFFFD; (*aktu&#xFFFD; (*aktu&#xFFFD; (*aktu&#xFFFD; (*aktu&#xFFFD; (*aktu&#xFFFD; (*aktu&#xFFFD; (*aktu&#xFFFD; (*aktu&#xFFFD; (*aktu&#xFFFD; (*aktu&#xFFFD; (*aktu&#xFFFD; (*aktu&#xFFFD; (*aktu&#xFFFD; (*aktu&#xFFFD; (*aktu&#xFFFD; (*aktu&#xFFFD; (*aktu&#xFFFD; (*aktu&#xFFFD; (*aktu&#xFFFD; (*aktu&#xFFFD; (*aktu&#xFFFD; (*aktu&#xFFFD; (*aktu&#xFFFD; (*aktu&#xFFFD; (*aktu&#xFFFD; (*aktu&#xFFFD; (*aktu&#xFFFD; (*aktu&#xFFFD; (*aktu&#xFFFD; (*aktu&#xFFFD; (*aktu&#xFFFD; (*aktu&#xFFFD; (*aktu&#xFFFD; (*aktu&#xFFFD; (*aktu&#xFFFD; (*aktu&#xFFFD; (*aktu&#xFFFD; (*aktu&#xFFFD; (*aktu&#xFFFD; (*aktu&#xFFFD; (*aktu&#xFFFD; (*aktu&#xFFFD; (*aktu&#xFFFD; (*aktu&#xFFFD; (*aktu&#xFFFD; (*aktu&#xFFFD; (*aktu&#xFFFD; (*aktu&#xFFFD; (*aktu&#xFFFD; (*aktu&#xFFFD; (*aktu&#xFFFD; (*aktu&#xFFFD; (*aktu&#xFFFD; (*aktu&#xFFFD; (*aktu&#xFFFD; (*aktu&#xFFFD; (*aktu&#xFFFD; (*aktu&#xFFFD; (*aktu&#xFFFD; (*aktu&#xFFFD; (*aktu&#xFFFD; (*aktu&#xFFFD; (*aktu&#xFFFD; (*aktu&#xFFFD; (*aktu&#xFFFD; (*aktu&#xFFFD; (*aktu&#xFFFD; (*aktu&#xFFFD; (*aktu&#xFFFD; (*aktu&#xFFFD; (*aktu&#xFFFD; (*aktu&#xFFFD; (*aktu&#xFFFD; (*aktu&#xFFFD; (*aktu&#xFFFD; (*aktu&#xFFFD; (*aktu&#xFFFD; (*aktu&#xFFFD; (*aktu&#xFFFD; (*aktu&#xFFFD; (*aktu&#xFFFD; (*aktu&#xFFFD; (*aktu&#xFFFD; (*aktu&#xFFFD; (*aktu&#xFFFD; (*aktu&#xFFFD; (*aktu&#xFFFD; (*aktu&#xFFFD; (*aktu&#xFFFD; (*aktu&#xFFFD; (*aktu&#xFFFD; (*aktu&#xFFFD; (*aktu&#xFFFD; (*aktu&#xFFFD; (*aktu&#xFFFD; (*aktu&#xFFFD; (*aktu&#xFFFD; (*aktu&#xFFFD; (*aktu&#xFFFD; (*aktu&#xFFFD; (*aktu&#xFFFD; (*aktu&#xFFFD; (*aktu&#xFFFD; (*aktu&#xFFFD; (*aktu&#xFFFD; (*aktu&#xFFFD; (*aktu&#xFFFD; (*aktu&#xFFFD; (*aktu&#xFFFD; (*aktu&#xFFFD; (*aktu&#xFFFD; (*aktu&#xFFFD; (*aktu&#xFFFD; (*aktu&#xFFFD; (*aktu&#xFFFD; (*aktu&#xFFFD; (*aktu&#xFFFD; (*aktu&#xFFFD; (*aktu&#xFFFD; (*aktu&#xFFFD; (*aktu&#xFFFD; (*aktu&#xFFFD; (*aktu&#xFFFD; (*aktu&#xFFFD; (*aktu&#xFFFD; (*aktu&#xFFFD; (*aktu&#xFFFD; (*aktu&#xFFFD; (*aktu&#xFFFD; (*aktu&#xFFFD; (*aktu&#xFFFD; (*aktu&#xFFFD; (*aktu&#xFFFD; (*aktu&#xFFFD; (*aktu&#xFFFD; (*aktu&#xFFFD; (*aktu&#xFFFD; (*aktu&#xFFFD; (*aktu&#xFFFD; (*aktu&#xFFFD; (*aktu&#xFFFD; (*aktu&#xFFFD; (*aktu&#xFFFD; (*aktu&#xFFFD; (*aktu&#xFFFD; (*aktu&#xFFFD; (*aktu&#xFFFD; (*aktu&#xFFFD; (*aktu&#xFFFD; (*aktu&#xFFFD; (*aktu&#xFFFD; (*aktu&#xFFFD; (*aktu&#xFFFD; (*aktu&#xFFFD; (*aktu&#xFFFD; (*aktu&#xFFFD; (*aktu&#xFFFD; (*aktu&#xFFFD; (*aktu&#xFFFD; (*aktu&#xFFFD; (*aktu&#xFFFD; (*aktu&#xFFFD; (*aktu&#xFFFD; (*aktu&#xFFFD; (*aktu&#xFFFD; (*aktu&#xFFFD; (*aktu&#xFFFD; (*aktu&#xFFFD; (*aktu&#xFFFD; (*aktu&#xFFFD; (*aktu&#xFFFD; (*aktu&#xFFFD; (*aktu&#xFFFD; (*aktu&#xFFFD; (*aktu&#xFFFD; (*aktu&#xFFFD; (*aktu&#xFFFD; (*aktu&#xFFFD; (*aktu&#xFFFD; (*aktu&#xFFFD; (*aktu&#xFFFD; (*aktu&#xFFFD; (*aktu&#xFFFD; (*aktu&#xFFFD; (*aktu&#xFFFD; (*aktu&#xFFFD; (*aktu&#xFFFD; (*aktu&#xFFFD; (*aktu&#xFFFD; (*aktu&#xFFFD; (*aktu&#xFFFD; (*aktu&#xFFFD; (*aktu&#xFFFD; (*aktu&#xFFFD; (*aktu&#xFFFD; (*aktu&#xFFFD; (*aktu&#xFFFD; (*aktu&#xFFFD; (*aktu&#xFFFD; (*aktu&#xFFFD; (*aktu&#xFFFD; (*aktu&#xFFFD; (*aktu&#xFFFD; (*aktu&#xFFFD; (*aktu&#xFFFD; (*aktu&#xFFFD; (*aktu&#xFFFD; (*aktu&#xFFFD; (*aktu&#xFFFD; (*aktu&#xFFFD; (*aktu&#xFFFD; (*aktu&#xFFFD; (*aktu&#xFFFD; (*aktu&#xFFFD; (*aktu&#xFFFD; (*aktu&#xFFFD; (*aktu&#xFFFD; (*aktu&#xFFFD; (*aktu&#xFFFD; (*aktu&#xFFFD; (*aktu&#xFFFD; (*aktu&#xFFFD; (*aktu&#xFFFD; (*aktu&#xFFFD; (*aktu&#xFFFD; (*aktu&#xFFFD; (*aktu&#xFFFD; (*aktu&#xFFFD; (*aktu&#xFFFD; (*aktu&#xFFFD; (*aktu&#xFFFD; (*aktu&#xFFFD; (*aktu&#xFFFD; (*aktu&#xFFFD; (*aktu&#xFFFD; (*aktu&#xFFFD; (*aktu&#xFFFD; (*aktu&#xFFFD; (*aktu&#xFFFD; (*aktu&#xFFFD; (*aktu&#xFFFD; (*aktu&#xFFFD; (*aktu&#xFFFD; (*aktu&#xFFFD; (*aktu&#xFFFD; (*aktu&#xFFFD; (*aktu&#xFFFD; (*aktu&#xFFFD; (*aktu&#xFFFD; (*aktu&#xFFFD; (*aktu&#xFFFD; (*aktu&#xFFFD; (*aktu&#xFFFD; (*aktu&#xFFFD; (*aktu&#xFFFD; (*aktu&#xFFFD; (*aktu&#xFFFD; (*aktu&#xFFFD; (*aktu&#xFFFD; (*aktu&#xFFFD; (*aktu&#xFFFD; (*aktu&#xFFFD; (*aktu&#xFFFD; (*aktu&#xFFFD; (*aktu&#xFFFD; (*aktu&#xFFFD; (*aktu&#xFFFD; (*aktu&#xFFFD; (*aktu&#xFFFD; (*aktu&#xFFFD; (*aktu&#xFFFD; (*aktu&#xFFFD; (*aktu&#xFFFD; (*aktu&#xFFFD; (*aktu&#xFFFD; (*aktu&#xFFFD; (*aktu&#xFFFD; (*aktu&#xFFFD; (*aktu&#xFFFD; (*aktu&#xFFFD; (*aktu&#xFFFD; (*aktu&#xFFFD; (*aktu&#xFFFD; (*aktu&#xFFFD; (*aktu&#xFFFD; (*aktu&#xFFFD; (*aktu&#xFFFD; (*aktu&#xFFFD; (*aktu&#xFFFD; (*aktu&#xFFFD; (*aktu&#xFFFD; (*aktu&#xFFFD; (*aktu&#xFFFD; (*aktu&#xFFFD; (*aktu&#xFFFD; (*aktu&#xFFFD; (*aktu&#xFFFD; (*aktu&#xFFFD; (*aktu&#xFFFD; (*aktu&#xFFFD; (*aktu&#xFFFD; (*aktu&#xFFFD; (*aktu&#xFFFD; (*aktu&#xFFFD; (*aktu&#xFFFD; (*aktu&#xFFFD; (*aktu&#xFFFD; (*aktu&#xFFFD; (*aktu&#xFFFD; (*aktu&#xFFFD; (*aktu&#xFFFD; (*aktu&#xFFFD; (*aktu&#xFFFD; (*aktu&#xFFFD; (*aktu&#xFFFD; (*aktu&#xFFFD; (*aktu&#xFFFD; (*aktu&#xFFFD; (*aktu&#xFFFD; (*aktu&#xFFFD; (*aktu&#xFFFD; (*aktu&#xFFFD; (*aktu&#xFFFD; (*aktu&#xFFFD; (*aktu&#xFFFD; (*aktu&#xFFFD; (*aktu&#xFFFD; (*aktu&#xFFFD; (*aktu&#xFFFD; (*aktu&#xFFFD; (*aktu&#xFFFD; (*aktu&#xFFFD; (*aktu&#xFFFD; (*aktu&#xFFFD; (*aktu&#xFFFD; (*aktu&#xFFFD; (*aktu&#xFFFD; (*aktu&#xFFFD; (*aktu&#xFFFD; (*aktu&#xFFFD; (*aktu&#xFFFD; (*aktu&#xFFFD; (*aktu&#xFFFD; (*aktu&#xFFFD; (*aktu&#xFFFD; (*aktu&#xFFFD; (*aktu&#xFFFD; (*aktu&#xFFFD; (*aktu&#xFFFD; (*aktu&#xFFFD; (*aktu&#xFFFD; (*aktu&#xFFFD; (*aktu&#xFFFD; (*aktu&#xFFFD; (*aktu&#xFFFD; (*aktu&#xFFFD; (*aktu&#xFFFD; (*aktu&#xFFFD; (*aktu&#xFFFD; (*aktu&#xFFFD; (*aktu&#xFFFD; (*aktu&#xFFFD; (*aktu&#xFFFD; (*aktu&#xFFFD; (*aktu&#xFFFD; (*aktu&#xFFFD; (*aktu&#xFFFD; (*aktu&#xFFFD; (*aktu&#xFFFD; (*aktu&#xFFFD; (*aktu&#xFFFD; (*aktu&#xFFFD; (*aktu&#xFFFD; (*aktu&#xFFFD; (*aktu&#xFFFD; (*aktu&#xFFFD; (*aktu&#xFFFD; (*aktu&#xFFFD; (*aktu&#xFFFD; (*aktu&#xFFFD; (*aktu&#xFFFD; (*aktu&#xFFFD; (*aktu&#xFFFD; (*aktu&#xFFFD; (*aktu&#xFFFD; (*aktu&#xFFFD; (*aktu&#xFFFD; (*aktu&#xFFFD; (*aktu&#xFFFD; (*aktu&#xFFFD; (*aktu&#xFFFD; (*aktu&#xFFFD; (*aktu&#xFFFD; (*aktu&#xFFFD; (*aktu&#xFFFD; (*aktu&#xFFFD; (*aktu&#xFFFD; (*aktu&#xFFFD; (*aktu&#xFFFD; (*aktu&#xFFFD; (*aktu&#xFFFD; (*aktu&#xFFFD; (*aktu&#xFFFD; (*aktu&#xFFFD; (*aktu&#xFFFD; (*aktu&#xFFFD; (*aktu&#xFFFD; (*aktu&#xFFFD; (*aktu&#xFFFD; (*aktu&#xFFFD; (*aktu&#xFFFD; (*aktu&#xFFFD; (*aktu&#xFFFD; (*aktu&#xFFFD; (*aktu&#xFFFD; (*aktu&#xFFFD; (*aktu&#xFFFD; (*aktu&#xFFFD; (*aktu&#xFFFD; (*aktu&#xFFFD; (*aktu&#xFFFD; (*aktu&#xFFFD; (*aktu&#xFFFD; (*aktu&#xFFFD; (*aktu&#xFFFD; (*aktu&#xFFFD; (*aktu&#xFFFD; (*aktu&#xFFFD; (*aktu&#xFFFD; (*aktu&#xFFFD; (*aktu&#xFFFD; (*aktu&#xFFFD; (*aktu&#xFFFD; (*aktu&#xFFFD; (*aktu&#xFFFD; (*aktu&#xFFFD; (*aktu&#xFFFD; (*aktu&#xFFFD; (*aktu&#xFFFD; (*aktu&#xFFFD; (*aktu&#xFFFD; (*aktu&#xFFFD; (*aktu&#xFFFD; (*aktu&#xFFFD; (*aktu&#xFFFD; (*aktu&#xFFFD; (*aktu&#xFFFD; (*aktu&#xFFFD; (*aktu&#xFFFD; (*aktu&#xFFFD; (*aktu&#xFFFD; (*aktu&#xFFFD; (*aktu&#xFFFD; (*aktu&#xFFFD; (*aktu&#xFFFD; (*aktu&#xFFFD; (*aktu&#xFFFD; (*aktu&#xFFFD; (*aktu&#xFFFD; (*aktu&#xFFFD; (*aktu&#xFFFD; (*aktu&#xFFFD; (*aktu&#xFFFD; (*aktu&#xFFFD; (*aktu&#xFFFD; (*aktu&#xFFFD; (*aktu&#xFFFD; (*aktu&#xFFFD; (*aktu&#xFFFD; (*aktu&#xFFFD; (*aktu&#xFFFD; (*aktu&#xFFFD; (*aktu&#xFFFD; (*aktu&#xFFFD; (*aktu&#xFFFD; (*aktu&#xFFFD; (*aktu&#xFFFD; (*aktu&#xFFFD; (*aktu&#xFFFD; (*aktu&#xFFFD; (*aktu&#xFFFD; (*aktu&#xFFFD; (*aktu&#xFFFD; (*aktu&#xFFFD; (*aktu&#xFFFD; (*aktu&#xFFFD; (*aktu&#xFFFD; (*aktu&#xFFFD; (*aktu&#xFFFD; (*aktu&#xFFFD; (*aktu&#xFFFD; (*aktu&#xFFFD; (*aktu&#xFFFD; (*aktu&#xFFFD; (*aktu&#xFFFD; (*aktu&#xFFFD; (*aktu&#xFFFD; (*aktu&#xFFFD; (*aktu&#xFFFD; (*aktu&#xFFFD; (*aktu&#xFFFD; (*aktu&#xFFFD; (*aktu&#xFFFD; (*aktu&#xFFFD; (*aktu&#xFFFD; (*aktu&#xFFFD; (*aktu&#xFFFD; (*aktu&#xFFFD; (*aktu&#xFFFD; (*aktu&#xFFFD; (*aktu&#xFFFD; (*aktu&#xFFFD; (*aktu&#xFFFD; (*aktu&#xFFFD; (*aktu&#xFFFD; (*aktu&#xFFFD; (*aktu&#xFFFD; (*aktu&#xFFFD; (*aktu&#xFFFD; (*aktu&#xFFFD; (*aktu&#xFFFD; (*aktu&#xFFFD; (*aktu&#xFFFD; (*aktu&#xFFFD; (*aktu&#xFFFD; (*aktu&#xFFFD; (*aktu&#xFFFD; (*aktu&#xFFFD; (*aktu&#xFFFD; (*aktu&#xFFFD; (*aktu&#xFFFD; (*aktu&#xFFFD; (*aktu&#xFFFD; (*aktu&#xFFFD; (*aktu&#xFFFD; (*aktu&#xFFFD; (*aktu&#xFFFD; (*aktu&#xFFFD; (*aktu&#xFFFD; (*aktu&#xFFFD; (*aktu&#xFFFD; (*aktu&#xFFFD; (*aktu&#xFFFD; (*aktu&#xFFFD; (*aktu&#xFFFD; (*aktu&#xFFFD; (*aktu&#xFFFD; (*aktu&#xFFFD; (*aktu&#xFFFD; (*aktu&#xFFFD; (*aktu&#xFFFD; (*aktu&#xFFFD; (*aktu&#xFFFD; (*aktu&#xFFFD; (*aktu&#xFFFD; (*aktu&#xFFFD; (*aktu&#xFFFD; (*aktu&#xFFFD; (*aktu&#xFFFD; (*aktu&#xFFFD; (*aktu&#xFFFD; (*aktu&#xFFFD; (*aktu&#xFFFD; (*aktu&#xFFFD; (*aktu&#xFFFD; (*aktu&#xFFFD; (*aktu&#xFFFD; (*aktu&#xFFFD; (*aktu&#xFFFD; (*aktu&#xFFFD; (*aktu&#xFFFD; (*aktu&#xFFFD; (*aktu&#xFFFD; (*aktu&#xFFFD; (*aktu&#xFFFD; (*aktu&#xFFFD; (*aktu&#xFFFD; (*aktu&#xFFFD; (*aktu&#xFFFD; (*aktu&#xFFFD; (*aktu&#xFFFD; (*aktu&#xFFFD; (*aktu&#xFFFD; (*aktu&#xFFFD; (*aktu&#xFFFD; (*aktu&#xFFFD; (*aktu&#xFFFD; (*aktu&#xFFFD; (*aktu&#xFFFD; (*aktu&#xFFFD; (*aktu&#xFFFD; (*aktu&#xFFFD; (*aktu&#xFFFD; (*aktu&#xFFFD; (*aktu&#xFFFD; (*aktu&#xFFFD; (*aktu&#xFFFD; (*aktu&#xFFFD; (*aktu&#xFFFD; (*aktu&#xFFFD; (*aktu&#xFFFD; (*aktu&#xFFFD; (*aktu&#xFFFD; (*aktu&#xFFFD; (*aktu&#xFFFD; (*aktu&#xFFFD; (*aktu&#xFFFD; (*aktu&#xFFFD; (*aktu&#xFFFD; (*aktu&#xFFFD; (*aktu&#xFFFD; (*aktu&#xFFFD; (*aktu&#xFFFD; (*aktu&#xFFFD; (*aktu&#xFFFD; (*aktu&#xFFFD; (*aktu&#xFFFD; (*aktu&#xFFFD; (*aktu&#xFFFD; (*aktu&#xFFFD; (*aktu&#xFFFD; (*aktu&#xFFFD; (*aktu&#xFFFD; (*aktu&#xFFFD; (*aktu&#xFFFD; (*aktu&#xFFFD; (*aktu&#xFFFD; (*aktu&#xFFFD; (*aktu&#xFFFD; (*aktu&#xFFFD; (*aktu&#xFFFD; (*aktu&#xFFFD; (*aktu&#xFFFD; (*aktu&#xFFFD; (*aktu&#xFFFD; (*aktu&#xFFFD; (*aktu&#xFFFD; (*aktu&#xFFFD; (*aktu&#xFFFD; (*aktu&#xFFFD; (*aktu&#xFFFD; (*aktu&#xFFFD; (*aktu&#xFFFD; (*aktu&#xFFFD; (*aktu&#xFFFD; (*aktu&#xFFFD; (*aktu&#xFFFD; (*aktu&#xFFFD; (*aktu&#xFFFD; (*aktu&#xFFFD; (*aktu&#xFFFD; (*aktu&#xFFFD; (*aktu&#xFFFD; (*aktu&#xFFFD; (*aktu&#xFFFD; (*aktu&#xFFFD; (*aktu&#xFFFD; (*aktu&#xFFFD; (*aktu&#xFFFD; (*aktu&#xFFFD; (*aktu&#xFFFD; (*aktu&#xFFFD; (*aktu&#xFFFD; (*aktu&#xFFFD; (*aktu&#xFFFD; (*aktu&#xFFFD; (*aktu&#xFFFD; (*aktu&#xFFFD; (*aktu&#xFFFD; (*aktu&#xFFFD; (*aktu&#xFFFD; (*aktu&#xFFFD; (*aktu&#xFFFD; (*aktu&#xFFFD; (*aktu&#xFFFD; (*aktu&#xFFFD; (*aktu&#xFFFD; (*aktu&#xFFFD; (*aktu&#xFFFD; (*aktu&#xFFFD; (*aktu&#xFFFD; (*aktu&#xFFFD; (*aktu&#xFFFD; (*aktu&#xFFFD; (*aktu&#xFFFD; (*aktu&#xFFFD; (*aktu&#xFFFD; (*aktu&#xFFFD; (*aktu&#xFFFD; (*aktu&#xFFFD; (*aktu&#xFFFD; (*aktu&#xFFFD; (*aktu&#xFFFD; (*aktu&#xFFFD; (*aktu&#xFFFD; (*aktu&#xFFFD; (*aktu&#xFFFD; (*aktu&#xFFFD; (*aktu&#xFFFD; (*aktu&#xFFFD; (*aktu&#xFFFD; (*aktu&#xFFFD; (*aktu&#xFFFD; (*aktu&#xFFFD; (*aktu&#xFFFD; (*aktu&#xFFFD; (*aktu&#xFFFD; (*aktu&#xFFFD; (*aktu&#xFFFD; (*aktu&#xFFFD; (*aktu&#xFFFD; (*aktu&#xFFFD; (*aktu&#xFFFD; (*aktu&#xFFFD; (*aktu&#xFFFD; (*aktu&#xFFFD; (*aktu&#xFFFD; (*aktu&#xFFFD; (*aktu&#xFFFD; (*aktu&#xFFFD; (*aktu&#xFFFD; (*aktu&#xFFFD; (*aktu&#xFFFD; (*aktu&#xFFFD; (*aktu&#xFFFD; (*aktu&#xFFFD; (*aktu&#xFFFD; (*aktu&#xFFFD; (*aktu&#xFFFD; (*aktu&#xFFFD; (*aktu&#xFFFD; (*aktu&#xFFFD; (*aktu&#xFFFD; (*aktu&#xFFFD; (*aktu&#xFFFD; (*aktu&#xFFFD; (*aktu&#xFFFD; (*aktu&#xFFFD; (*aktu&#xFFFD; (*aktu&#xFFFD; (*aktu&#xFFFD; (*aktu&#xFFFD; (*aktu&#xFFFD; (*aktu&#xFFFD; (*aktu&#xFFFD; (*aktu&#xFFFD; (*aktu&#xFFFD; (*aktu&#xFFFD; (*aktu&#xFFFD; (*aktu&#xFFFD; (*aktu&#xFFFD; (*aktu&#xFFFD; (*aktu&#xFFFD; (*aktu&#xFFFD; (*aktu&#xFFFD; (*aktu&#xFFFD; (*aktu&#xFFFD; (*aktu&#xFFFD; (*aktu&#xFFFD; (*aktu&#xFFFD; (*aktu&#xFFFD; (*aktu&#xFFFD; (*aktu&#xFFFD; (*aktu&#xFFFD; (*aktu&#xFFFD; (*aktu&#xFFFD; (*aktu&#xFFFD; (*aktu&#xFFFD; (*aktu&#xFFFD; (*aktu&#xFFFD; (*aktu&#xFFFD; (*aktu&#xFFFD; (*aktu&#xFFFD; (*aktu&#xFFFD; (*aktu&#xFFFD; (*aktu&#xFFFD; (*aktu&#xFFFD; (*aktu&#xFFFD; (*aktu&#xFFFD; (*aktu&#xFFFD; (*aktu&#xFFFD; (*aktu&#xFFFD; (*aktu&#xFFFD; (*aktu&#xFFFD; (*aktu&#xFFFD; (*aktu&#xFFFD; (*aktu&#xFFFD; (*aktu&#xFFFD; (*aktu&#xFFFD; (*aktu&#xFFFD; (*aktu&#xFFFD; (*aktu&#xFFFD; (*aktu&#xFFFD; (*aktu&#xFFFD; (*aktu&#xFFFD; (*aktu&#xFFFD; (*aktu&#xFFFD; (*aktu&#xFFFD; (*aktu&#xFFFD; (*aktu&#xFFFD; (*aktu&#xFFFD; (*aktu&#xFFFD; (*aktu&#xFFFD; (*aktu&#xFFFD; (*aktu&#xFFFD; (*aktu&#xFFFD; (*aktu&#xFFFD; (*aktu&#xFFFD; (*aktu&#xFFFD; (*aktu&#xFFFD; (*aktu&#xFFFD; (*aktu&#xFFFD; (*aktu&#xFFFD; (*aktu&#xFFFD; (*aktu&#xFFFD; (*aktu&#xFFFD; (*aktu&#xFFFD; (*aktu&#xFFFD; (*aktu&#xFFFD; (*aktu&#xFFFD; (*aktu&#xFFFD; (*aktu&#xFFFD; (*aktu&#xFFFD; (*aktu&#xFFFD; (*aktu&#xFFFD; (*aktu&#xFFFD; (*aktu&#xFFFD; (*aktu&#xFFFD; (*aktu&#xFFFD; (*aktu&#xFFFD; (*aktu&#xFFFD; (*aktu&#xFFFD; (*aktu&#xFFFD; (*aktu&#xFFFD; (*aktu&#xFFFD; (*aktu&#xFFFD; (*aktu&#xFFFD; (*aktu&#xFFFD; (*aktu&#xFFFD; (*aktu&#xFFFD; (*aktu&#xFFFD; (*aktu&#xFFFD; (*aktu&#xFFFD; (*aktu&#xFFFD; (*aktu&#xFFFD; (*aktu&#xFFFD; (*aktu&#xFFFD; (*aktu&#xFFFD; (*aktu&#xFFFD; (*aktu&#xFFFD; (*aktu&#xFFFD; (*aktu&#xFFFD; (*aktu&#xFFFD; (*aktu&#xFFFD; (*aktu&#xFFFD; (*aktu&#xFFFD; (*aktu&#xFFFD; (*aktu&#xFFFD; (*aktu&#xFFFD; (*aktu&#xFFFD; (*aktu&#xFFFD; (*aktu&#xFFFD; (*aktu&#xFFFD; (*aktu&#xFFFD; (*aktu&#xFFFD; (*aktu&#xFFFD; (*aktu&#xFFFD; (*aktu&#xFFFD; (*aktu&#xFFFD; (*aktu&#xFFFD; (*aktu&#xFFFD; (*aktu&#xFFFD; (*aktu&#xFFFD; (*aktu&#xFFFD; (*aktu&#xFFFD; (*aktu&#xFFFD; (*aktu&#xFFFD; (*aktu&#xFFFD; (*aktu&#xFFFD; (*aktu&#xFFFD; (*aktu&#xFFFD; (*aktu&#xFFFD; (*aktu&#xFFFD; (*aktu&#xFFFD; (*aktu&#xFFFD; (*aktu&#xFFFD; (*aktu&#xFFFD; (*aktu&#xFFFD; (*aktu&#xFFFD; (*aktu&#xFFFD; (*aktu&#xFFFD; (*aktu&#xFFFD; (*aktu&#xFFFD; (*aktu&#xFFFD; (*aktu&#xFFFD; (*aktu&#xFFFD; (*aktu&#xFFFD; (*aktu&#xFFFD; (*aktu&#xFFFD; (*aktu&#xFFFD; (*aktu&#xFFFD; (*aktu&#xFFFD; (*aktu&#xFFFD; (*aktu&#xFFFD; (*aktu&#xFFFD; (*aktu&#xFFFD; (*aktu&#xFFFD; (*aktu&#xFFFD; (*aktu&#xFFFD; (*aktu&#xFFFD; (*aktu&#xFFFD; (*aktu&#xFFFD; (*aktu&#xFFFD; (*aktu&#xFFFD; (*aktu&#xFFFD; (*aktu&#xFFFD; (*aktu&#xFFFD; (*aktu&#xFFFD; (*aktu&#xFFFD; (*aktu&#xFFFD; (*aktu&#xFFFD; (*aktu&#xFFFD; (*aktu&#xFFFD; (*aktu&#xFFFD; (*aktu&#xFFFD; (*aktu&#xFFFD; (*aktu&#xFFFD; (*aktu&#xFFFD; (*aktu&#xFFFD; (*aktu&#xFFFD; (*aktu&#xFFFD; (*aktu&#xFFFD; (*aktu&#xFFFD; (*aktu&#xFFFD; (*aktu&#xFFFD; (*aktu&#xFFFD; (*aktu&#xFFFD; (*aktu&#xFFFD; (*aktu&#xFFFD; (*aktu&#xFFFD; (*aktu&#xFFFD; (*aktu&#xFFFD; (*aktu&#xFFFD; (*aktu&#xFFFD; (*aktu&#xFFFD; (*aktu&#xFFFD; (*aktu&#xFFFD; (*aktu&#xFFFD; (*aktu&#xFFFD; (*aktu&#xFFFD; (*aktu&#xFFFD; (*aktu&#xFFFD; (*aktu&#xFFFD; (*aktu&#xFFFD; (*aktu&#xFFFD; (*aktu&#xFFFD; (*aktu&#xFFFD; (*aktu&#xFFFD; (*aktu&#xFFFD; (*aktu&#xFFFD; (*aktu&#xFFFD; (*aktu&#xFFFD; (*aktu&#xFFFD; (*aktu&#xFFFD; (*aktu&#xFFFD; (*aktu&#xFFFD; (*aktu&#xFFFD; (*aktu&#xFFFD; (*aktu&#xFFFD; (*aktu&#xFFFD; (*aktu&#xFFFD; (*aktu&#xFFFD; (*aktu&#xFFFD; (*aktu&#xFFFD; (*aktu&#xFFFD; (*aktu&#xFFFD; (*aktu&#xFFFD; (*aktu&#xFFFD; (*aktu&#xFFFD; (*aktu&#xFFFD; (*aktu&#xFFFD; (*aktu&#xFFFD; (*aktu&#xFFFD; (*aktu&#xFFFD; (*aktu&#xFFFD; (*aktu&#xFFFD; (*aktu&#xFFFD; (*aktu&#xFFFD; (*aktu&#xFFFD; (*aktu&#xFFFD; (*aktu&#xFFFD; (*aktu&#xFFFD; (*aktu&#xFFFD; (*aktu&#xFFFD; (*aktu&#xFFFD; (*aktu&#xFFFD; (*aktu&#xFFFD; (*aktu&#xFFFD; (*aktu&#xFFFD; (*aktu&#xFFFD; (*aktu&#xFFFD; (*aktu&#xFFFD; (*aktu&#xFFFD; (*aktu&#xFFFD; (*aktu&#xFFFD; (*aktu&#xFFFD; (*aktu&#xFFFD; (*aktu&#xFFFD; (*aktu&#xFFFD; (*aktu&#xFFFD; (*aktu&#xFFFD; (*aktu&#xFFFD; (*aktu&#xFFFD; (*aktu&#xFFFD; (*aktu&#xFFFD; (*aktu&#xFFFD; (*aktu&#xFFFD; (*aktu&#xFFFD; (*aktu&#xFFFD; (*aktu&#xFFFD; (*aktu&#xFFFD; (*aktu&#xFFFD; (*aktu&#xFFFD; (*aktu&#xFFFD; (*aktu&#xFFFD; (*aktu&#xFFFD; (*aktu&#xFFFD; (*aktu&#xFFFD; (*aktu&#xFFFD; (*aktu&#xFFFD; (*aktu&#xFFFD; (*aktu&#xFFFD; (*aktu&#xFFFD; (*aktu&#xFFFD; (*aktu&#xFFFD; (*aktu&#xFFFD; (*aktu&#xFFFD; (*aktu&#xFFFD; (*aktu&#xFFFD; (*aktu&#xFFFD; (*aktu&#xFFFD; (*aktu&#xFFFD; (*aktu&#xFFFD; (*aktu&#xFFFD; (*aktu&#xFFFD; (*aktu&#xFFFD; (*aktu&#xFFFD; (*aktu&#xFFFD; (*aktu&#xFFFD; (*aktu&#xFFFD; (*aktu&#xFFFD; (*aktu&#xFFFD; (*aktu&#xFFFD; (*aktu&#xFFFD; (*aktu&#xFFFD; (*aktu&#xFFFD; (*aktu&#xFFFD; (*aktu&#xFFFD; (*aktu&#xFFFD; (*aktu&#xFFFD; (*aktu&#xFFFD; (*aktu&#xFFFD; (*aktu&#xFFFD; (*aktu&#xFFFD; (*aktu&#xFFFD; (*aktu&#xFFFD; (*aktu&#xFFFD; (*aktu&#xFFFD; (*aktu&#xFFFD; (*aktu&#xFFFD; (*aktu&#xFFFD; (*aktu&#xFFFD; (*aktu&#xFFFD; (*aktu&#xFFFD; (*aktu&#xFFFD; (*aktu&#xFFFD; (*aktu&#xFFFD; (*aktu&#xFFFD; (*aktu&#xFFFD; (*aktu&#xFFFD; (*aktu&#xFFFD; (*aktu&#xFFFD; (*aktu&#xFFFD; (*aktu&#xFFFD; (*aktu&#xFFFD; (*aktu&#xFFFD; (*aktu&#xFFFD; (*aktu&#xFFFD; (*aktu&#xFFFD; (*aktu&#xFFFD; (*aktu&#xFFFD; (*aktu&#xFFFD; (*aktu&#xFFFD; (*aktu&#xFFFD; (*aktu&#xFFFD; (*aktu&#xFFFD; (*aktu&#xFFFD; (*aktu&#xFFFD; (*aktu&#xFFFD; (*aktu&#xFFFD; (*aktu&#xFFFD; (*aktu&#xFFFD; (*aktu&#xFFFD; (*aktu&#xFFFD; (*aktu&#xFFFD; (*aktu&#xFFFD; (*aktu&#xFFFD; (*aktu&#xFFFD; (*aktu&#xFFFD; (*aktu&#xFFFD; (*aktu&#xFFFD; (*aktu&#xFFFD; (*aktu&#xFFFD; (*aktu&#xFFFD; (*aktu&#xFFFD; (*aktu&#xFFFD; (*aktu&#xFFFD; (*aktu&#xFFFD; (*aktu&#xFFFD; (*aktu&#xFFFD; (*aktu&#xFFFD; (*aktu&#xFFFD; (*aktu&#xFFFD; (*aktu&#xFFFD; (*aktu&#xFFFD; (*aktu&#xFFFD; (*aktu&#xFFFD; (*aktu&#xFFFD; (*aktu&#xFFFD; (*aktu&#xFFFD; (*aktu&#xFFFD; (*aktu&#xFFFD; (*aktu&#xFFFD; (*aktu&#xFFFD; (*aktu&#xFFFD; (*aktu&#xFFFD; (*aktu&#xFFFD; (*aktu&#xFFFD; (*aktu&#xFFFD; (*aktu&#xFFFD; (*aktu&#xFFFD; (*aktu&#xFFFD; (*aktu&#xFFFD; (*aktu&#xFFFD; (*aktu&#xFFFD; (*aktu&#xFFFD; (*aktu&#xFFFD; (*aktu&#xFFFD; (*aktu&#xFFFD; (*aktu&#xFFFD; (*aktu&#xFFFD; (*aktu&#xFFFD; (*aktu&#xFFFD; (*aktu&#xFFFD; (*aktu&#xFFFD; (*aktu&#xFFFD; (*aktu&#xFFFD; (*aktu&#xFFFD; (*aktu&#xFFFD; (*aktu&#xFFFD; (*aktu&#xFFFD; (*aktu&#xFFFD; (*aktu&#xFFFD; (*aktu&#xFFFD; (*aktu&#xFFFD; (*aktu&#xFFFD; (*aktu&#xFFFD; (*aktu&#xFFFD; (*aktu&#xFFFD; (*aktu&#xFFFD; (*aktu&#xFFFD; (*aktu&#xFFFD; (*aktu&#xFFFD; (*aktu&#xFFFD; (*aktu&#xFFFD; (*aktu&#xFFFD; (*aktu&#xFFFD; (*aktu&#xFFFD; (*aktu&#xFFFD; (*aktu&#xFFFD; (*aktu&#xFFFD; (*aktu&#xFFFD; (*aktu&#xFFFD; (*aktu&#xFFFD; (*aktu&#xFFFD; (*aktu&#xFFFD; (*aktu&#xFFFD; (*aktu&#xFFFD; (*aktu&#xFFFD; (*aktu&#xFFFD; (*aktu&#xFFFD; (*aktu&#xFFFD; (*aktu&#xFFFD; (*aktu&#xFFFD; (*aktu&#xFFFD; (*aktu&#xFFFD; (*aktu&#xFFFD; (*aktu&#xFFFD; (*aktu&#xFFFD; (*aktu&#xFFFD; (*aktu&#xFFFD; (*aktu&#xFFFD; (*aktu&#xFFFD; (*aktu&#xFFFD; (*aktu&#xFFFD; (*aktu&#xFFFD; (*aktu&#xFFFD; (*aktu&#xFFFD; (*aktu&#xFFFD; (*aktu&#xFFFD; (*aktu&#xFFFD; (*aktu&#xFFFD; (*aktu&#xFFFD; (*aktu&#xFFFD; (*aktu&#xFFFD; (*aktu&#xFFFD; (*aktu&#xFFFD; (*aktu&#xFFFD; (*aktu&#xFFFD; (*aktu&#xFFFD; (*aktu&#xFFFD; (*aktu&#xFFFD; (*aktu&#xFFFD; (*aktu&#xFFFD; (*aktu&#xFFFD; (*aktu&#xFFFD; (*aktu&#xFFFD; (*aktu&#xFFFD; (*aktu&#xFFFD; (*aktu&#xFFFD; (*aktu&#xFFFD; (*aktu&#xFFFD; (*aktu&#xFFFD; (*aktu&#xFFFD; (*aktu&#xFFFD; (*aktu&#xFFFD; (*aktu&#xFFFD; (*aktu&#xFFFD; (*aktu&#xFFFD; (*aktu&#xFFFD; (*aktu&#xFFFD; (*aktu&#xFFFD; (*aktu&#xFFFD; (*aktu&#xFFFD; (*aktu&#xFFFD; (*aktu&#xFFFD; (*aktu&#xFFFD; (*aktu&#xFFFD; (*aktu&#xFFFD; (*aktu&#xFFFD; (*aktu&#xFFFD; (*aktu&#xFFFD; (*aktu&#xFFFD; (*aktu&#xFFFD; (*aktu&#xFFFD; (*aktu&#xFFFD; (*aktu&#xFFFD; (*aktu&#xFFFD; (*aktu&#xFFFD; (*aktu&#xFFFD; (*aktu&#xFFFD; (*aktu&#xFFFD; (*aktu&#xFFFD; (*aktu&#xFFFD; (*aktu&#xFFFD; (*aktu&#xFFFD; (*aktu&#xFFFD; (*aktu&#xFFFD; (*aktu&#xFFFD; (*aktu&#xFFFD; (*aktu&#xFFFD; (*aktu&#xFFFD; (*aktu&#xFFFD; (*aktu&#xFFFD; (*aktu&#xFFFD; (*aktu&#xFFFD; (*aktu&#xFFFD; (*aktu&#xFFFD; (*aktu&#xFFFD; (*aktu&#xFFFD; (*aktu&#xFFFD; (*aktu&#xFFFD; (*aktu&#xFFFD; (*aktu&#xFFFD; (*aktu&#xFFFD; (*aktu&#xFFFD; (*aktu&#xFFFD; (*aktu&#xFFFD; (*aktu&#xFFFD; (*aktu&#xFFFD; (*aktu&#xFFFD; (*aktu&#xFFFD; (*aktu&#xFFFD; (*aktu&#xFFFD; (*aktu&#xFFFD; (*aktu&#xFFFD; (*aktu&#xFFFD; (*aktu&#xFFFD; (*aktu&#xFFFD; (*aktu&#xFFFD; (*aktu&#xFFFD; (*aktu&#xFFFD; (*aktu&#xFFFD; (*aktu&#xFFFD; (*aktu&#xFFFD; (*aktu&#xFFFD; (*aktu&#xFFFD; (*aktu&#xFFFD; (*aktu&#xFFFD; (*aktu&#xFFFD; (*aktu&#xFFFD; (*aktu&#xFFFD; (*aktu&#xFFFD; (*aktu&#xFFFD; (*aktu&#xFFFD; (*aktu&#xFFFD; (*aktu&#xFFFD; (*aktu&#xFFFD; (*aktu&#xFFFD; (*aktu&#xFFFD; (*aktu&#xFFFD; (*aktu&#xFFFD; (*aktu&#xFFFD; (*aktu&#xFFFD; (*aktu&#xFFFD; (*aktu&#xFFFD; (*aktu&#xFFFD; (*aktu&#xFFFD; (*aktu&#xFFFD; (*aktu&#xFFFD; (*aktu&#xFFFD; (*aktu&#xFFFD; (*aktu&#xFFFD; (*aktu&#xFFFD; (*aktu&#xFFFD; (*aktu&#xFFFD; (*aktu&#xFFFD; (*aktu&#xFFFD; (*aktu&#xFFFD; (*aktu&#xFFFD; (*aktu&#xFFFD; (*aktu&#xFFFD; (*aktu&#xFFFD; (*aktu&#xFFFD; (*aktu&#xFFFD; (*aktu&#xFFFD; (*aktu&#xFFFD; (*aktu&#xFFFD; (*aktu&#xFFFD; (*aktu&#xFFFD; (*aktu&#xFFFD; (*aktu&#xFFFD; (*aktu&#xFFFD; (*aktu&#xFFFD; (*aktu&#xFFFD; (*aktu&#xFFFD; (*aktu&#xFFFD; (*aktu&#xFFFD; (*aktu&#xFFFD; (*aktu&#xFFFD; (*aktu&#xFFFD; (*aktu&#xFFFD; (*aktu&#xFFFD; (*aktu&#xFFFD; (*aktu&#xFFFD; (*aktu&#xFFFD; (*aktu&#xFFFD; (*aktu&#xFFFD; (*aktu&#xFFFD; (*aktu&#xFFFD; (*aktu&#xFFFD; (*aktu&#xFFFD; (*aktu&#xFFFD; (*aktu&#xFFFD; (*aktu&#xFFFD; (*aktu&#xFFFD; (*aktu&#xFFFD; (*aktu&#xFFFD; (*aktu&#xFFFD; (*aktu&#xFFFD; (*aktu&#xFFFD; (*aktu&#xFFFD; (*aktu&#xFFFD; (*aktu&#xFFFD; (*aktu&#xFFFD; (*aktu&#xFFFD; (*aktu&#xFFFD; (*aktu&#xFFFD; (*aktu&#xFFFD; (*aktu&#xFFFD; (*aktu&#xFFFD; (*aktu&#xFFFD; (*aktu&#xFFFD; (*aktu&#xFFFD; (*aktu&#xFFFD; (*aktu&#xFFFD; (*aktu&#xFFFD; (*aktu&#xFFFD; (*aktu&#xFFFD; (*aktu&#xFFFD; (*aktu&#xFFFD; (*aktu&#xFFFD; (*aktu&#xFFFD; (*aktu&#xFFFD; (*aktu&#xFFFD; (*aktu&#xFFFD; (*aktu&#xFFFD; (*aktu&#xFFFD; (*aktu&#xFFFD; (*aktu&#xFFFD; (*aktu&#xFFFD; (*aktu&#xFFFD; (*aktu&#xFFFD; (*aktu&#xFFFD; (*aktu&#xFFFD; (*aktu&#xFFFD; (*aktu&#xFFFD; (*aktu&#xFFFD; (*aktu&#xFFFD; (*aktu&#xFFFD; (*aktu&#xFFFD; (*aktu&#xFFFD; (*aktu&#xFFFD; (*aktu&#xFFFD; (*aktu&#xFFFD; (*aktu&#xFFFD; (*aktu&#xFFFD; (*aktu&#xFFFD; (*aktu&#xFFFD; (*aktu&#xFFFD; (*aktu&#xFFFD; (*aktu&#xFFFD; (*aktu&#xFFFD; (*aktu&#xFFFD; (*aktu&#xFFFD; (*aktu&#xFFFD; (*aktu&#xFFFD; (*aktu&#xFFFD; (*aktu&#xFFFD; (*aktu&#xFFFD; (*aktu&#xFFFD; (*aktu&#xFFFD; (*aktu&#xFFFD; (*aktu&#xFFFD; (*aktu&#xFFFD; (*aktu&#xFFFD; (*aktu&#xFFFD; (*aktu&#xFFFD; (*aktu&#xFFFD; (*aktu&#xFFFD; (*aktu&#xFFFD; (*aktu&#xFFFD; (*aktu&#xFFFD; (*aktu&#xFFFD; (*aktu&#xFFFD; (*aktu&#xFFFD; (*aktu&#xFFFD; (*aktu&#xFFFD; (*aktu&#xFFFD; (*aktu&#xFFFD; (*aktu&#xFFFD; (*aktu&#xFFFD; (*aktu&#xFFFD; (*aktu&#xFFFD; (*aktu&#xFFFD; (*aktu&#xFFFD; (*aktu&#xFFFD; (*aktu&#xFFFD; (*aktu&#xFFFD; (*aktu&#xFFFD; (*aktu&#xFFFD; (*aktu&#xFFFD; (*aktu&#xFFFD; (*aktu&#xFFFD; (*aktu&#xFFFD; (*aktu&#xFFFD; (*aktu&#xFFFD; (*aktu&#xFFFD; (*aktu&#xFFFD; (*aktu&#xFFFD; (*aktu&#xFFFD; (*aktu&#xFFFD; (*aktu&#xFFFD; (*aktu&#xFFFD; (*aktu&#xFFFD; (*aktu&#xFFFD; (*aktu&#xFFFD; (*aktu&#xFFFD; (*aktu&#xFFFD; (*aktu&#xFFFD; (*aktu&#xFFFD; (*aktu&#xFFFD; (*aktu&#xFFFD; (*aktu&#xFFFD; (*aktu&#xFFFD; (*aktu&#xFFFD; (*aktu&#xFFFD; (*aktu&#xFFFD; (*aktu&#xFFFD; (*aktu&#xFFFD; (*aktu&#xFFFD; (*aktu&#xFFFD; (*aktu&#xFFFD; (*aktu&#xFFFD; (*aktu&#xFFFD; (*aktu&#xFFFD; (*aktu&#xFFFD; (*aktu&#xFFFD; (*aktu&#xFFFD; (*aktu&#xFFFD; (*aktu&#xFFFD; (*aktu&#xFFFD; (*aktu&#xFFFD; (*aktu&#xFFFD; (*aktu&#xFFFD; (*aktu&#xFFFD; (*aktu&#xFFFD; (*aktu&#xFFFD; (*aktu&#xFFFD; (*aktu&#xFFFD; (*aktu&#xFFFD; (*aktu&#xFFFD; (*aktu&#xFFFD; (*aktu&#xFFFD; (*aktu&#xFFFD; (*aktu&#xFFFD; (*aktu&#xFFFD; (*aktu&#xFFFD; (*aktu&#xFFFD; (*aktu&#xFFFD; (*aktu&#xFFFD; (*aktu&#xFFFD; (*aktu&#xFFFD; (*aktu&#xFFFD; (*aktu&#xFFFD; (*aktu&#xFFFD; (*aktu&#xFFFD; (*aktu&#xFFFD; (*aktu&#xFFFD; (*aktu&#xFFFD; (*aktu&#xFFFD; (*aktu&#xFFFD; (*aktu&#xFFFD; (*aktu&#xFFFD; (*aktu&#xFFFD; (*aktu&#xFFFD; (*aktu&#xFFFD; (*aktu&#xFFFD; (*aktu&#xFFFD; (*aktu&#xFFFD; (*aktu&#xFFFD; (*aktu&#xFFFD; (*aktu&#xFFFD; (*aktu&#xFFFD; (*aktu&#xFFFD; (*aktu&#xFFFD; (*aktu&#xFFFD; (*aktu&#xFFFD; (*aktu&#xFFFD; (*aktu&#xFFFD; (*aktu&#xFFFD; (*aktu&#xFFFD; (*aktu&#xFFFD; (*aktu&#xFFFD; (*aktu&#xFFFD; (*aktu&#xFFFD; (*aktu&#xFFFD; (*aktu&#xFFFD; (*aktu&#xFFFD; (*aktu&#xFFFD; (*aktu&#xFFFD; (*aktu&#xFFFD; (*aktu&#xFFFD; (*aktu&#xFFFD; (*aktu&#xFFFD; (*aktu&#xFFFD; (*aktu&#xFFFD; (*aktu&#xFFFD; (*aktu&#xFFFD; (*aktu&#xFFFD; (*aktu&#xFFFD; (*aktu&#xFFFD; (*aktu&#xFFFD; (*aktu&#xFFFD; (*aktu&#xFFFD; (*aktu&#xFFFD; (*aktu&#xFFFD; (*aktu&#xFFFD; (*aktu&#xFFFD; (*aktu&#xFFFD; (*aktu&#xFFFD; (*aktu&#xFFFD; (*aktu&#xFFFD; (*aktu&#xFFFD; (*aktu&#xFFFD; (*aktu&#xFFFD; (*aktu&#xFFFD; (*aktu&#xFFFD; (*aktu&#xFFFD; (*aktu&#xFFFD; (*aktu&#xFFFD; (*aktu&#xFFFD; (*aktu&#xFFFD; (*aktu&#xFFFD; (*aktu&#xFFFD; (*aktu&#xFFFD; (*aktu&#xFFFD; (*aktu&#xFFFD; (*aktu&#xFFFD; (*aktu&#xFFFD; (*aktu&#xFFFD; (*aktu&#xFFFD; (*aktu&#xFFFD; (*aktu&#xFFFD; (*aktu&#xFFFD; (*aktu&#xFFFD; (*aktu&#xFFFD; (*aktu&#xFFFD; (*aktu&#xFFFD; (*aktu&#xFFFD; (*aktu&#xFFFD; (*aktu&#xFFFD; (*aktu&#xFFFD; (*aktu&#xFFFD; (*aktu&#xFFFD; (*aktu&#xFFFD; (*aktu&#xFFFD; (*aktu&#xFFFD; (*aktu&#xFFFD; (*aktu&#xFFFD; (*aktu&#xFFFD; (*aktu&#xFFFD; (*aktu&#xFFFD; (*aktu&#xFFFD; (*aktu&#xFFFD; (*aktu&#xFFFD; (*aktu&#xFFFD; (*aktu&#xFFFD; (*aktu&#xFFFD; (*aktu&#xFFFD; (*aktu&#xFFFD; (*aktu&#xFFFD; (*aktu&#xFFFD; (*aktu&#xFFFD; (*aktu&#xFFFD; (*aktu&#xFFFD; (*aktu&#xFFFD; (*aktu&#xFFFD; (*aktu&#xFFFD; (*aktu&#xFFFD; (*aktu&#xFFFD; (*aktu&#xFFFD; (*aktu&#xFFFD; (*aktu&#xFFFD; (*aktu&#xFFFD; (*aktu&#xFFFD; (*aktu&#xFFFD; (*aktu&#xFFFD; (*aktu&#xFFFD; (*aktu&#xFFFD; (*aktu&#xFFFD; (*aktu&#xFFFD; (*aktu&#xFFFD; (*aktu&#xFFFD; (*aktu&#xFFFD; (*aktu&#xFFFD; (*aktu&#xFFFD; (*aktu&#xFFFD; (*aktu&#xFFFD; (*aktu&#xFFFD; (*aktu&#xFFFD; (*aktu&#xFFFD; (*aktu&#xFFFD; (*aktu&#xFFFD; (*aktu&#xFFFD; (*aktu&#xFFFD; (*aktu&#xFFFD; (*aktu&#xFFFD; (*aktu&#xFFFD; (*aktu&#xFFFD; (*aktu&#xFFFD; (*aktu&#xFFFD; (*aktu&#xFFFD; (*aktu&#xFFFD; (*aktu&#xFFFD; (*aktu&#xFFFD; (*aktu&#xFFFD; (*aktu&#xFFFD; (*aktu&#xFFFD; (*aktu&#xFFFD; (*aktu&#xFFFD; (*aktu&#xFFFD; (*aktu&#xFFFD; (*aktu&#xFFFD; (*aktu&#xFFFD; (*aktu&#xFFFD; (*aktu&#xFFFD; (*aktu&#xFFFD; (*aktu&#xFFFD; (*aktu&#xFFFD; (*aktu&#xFFFD; (*aktu&#xFFFD; (*aktu&#xFFFD; (*aktu&#xFFFD; (*aktu&#xFFFD; (*aktu&#xFFFD; (*aktu&#xFFFD; (*aktu&#xFFFD; (*aktu&#xFFFD; (*aktu&#xFFFD; (*aktu&#xFFFD; (*aktu&#xFFFD; (*aktu&#xFFFD; (*aktu&#xFFFD; (*aktu&#xFFFD; (*aktu&#xFFFD; (*aktu&#xFFFD; (*aktu&#xFFFD; (*aktu&#xFFFD; (*aktu&#xFFFD; (*aktu&#xFFFD; (*aktu&#xFFFD; (*aktu&#xFFFD; (*aktu&#xFFFD; (*aktu&#xFFFD; (*aktu&#xFFFD; (*aktu&#xFFFD; (*aktu&#xFFFD; (*aktu&#xFFFD; (*aktu&#xFFFD; (*aktu&#xFFFD; (*aktu&#xFFFD; (*aktu&#xFFFD; (*aktu&#xFFFD; (*aktu&#xFFFD; (*aktu&#xFFFD; (*aktu&#xFFFD; (*aktu&#xFFFD; (*aktu&#xFFFD; (*aktu&#xFFFD; (*aktu&#xFFFD; (*aktu&#xFFFD; (*aktu&#xFFFD; (*aktu&#xFFFD; (*aktu&#xFFFD; (*aktu&#xFFFD; (*aktu&#xFFFD; (*aktu&#xFFFD; (*aktu&#xFFFD; (*aktu&#xFFFD; (*aktu&#xFFFD; (*aktu&#xFFFD; (*aktu&#xFFFD; (*aktu&#xFFFD; (*aktu&#xFFFD; (*aktu&#xFFFD; (*aktu&#xFFFD; (*aktu&#xFFFD; (*aktu&#xFFFD; (*aktu&#xFFFD; (*aktu&#xFFFD; (*aktu&#xFFFD; (*aktu&#xFFFD; (*aktu&#xFFFD; (*aktu&#xFFFD; (*aktu&#xFFFD; (*aktu&#xFFFD; (*aktu&#xFFFD; (*aktu&#xFFFD; (*aktu&#xFFFD; (*aktu&#xFFFD; (*aktu&#xFFFD; (*aktu&#xFFFD; (*aktu&#xFFFD; (*aktu&#xFFFD; (*aktu&#xFFFD; (*aktu&#xFFFD; (*aktu&#xFFFD; (*aktu&#xFFFD; (*aktu&#xFFFD; (*aktu&#xFFFD; (*aktu&#xFFFD; (*aktu&#xFFFD; (*aktu&#xFFFD; (*aktu&#xFFFD; (*aktu&#xFFFD; (*aktu&#xFFFD; (*aktu&#xFFFD; (*aktu&#xFFFD; (*aktu&#xFFFD; (*aktu&#xFFFD; (*aktu&#xFFFD; (*aktu&#xFFFD; (*aktu&#xFFFD; (*aktu&#xFFFD; (*aktu&#xFFFD; (*aktu&#xFFFD; (*aktu&#xFFFD; (*aktu&#xFFFD; (*aktu&#xFFFD; (*aktu&#xFFFD; (*aktu&#xFFFD; (*aktu&#xFFFD; (*aktu&#xFFFD; (*aktu&#xFFFD; (*aktu&#xFFFD; (*aktu&#xFFFD; (*aktu&#xFFFD; (*aktu&#xFFFD; (*aktu&#xFFFD; (*aktu&#xFFFD; (*aktu&#xFFFD; (*aktu&#xFFFD; (*aktu&#xFFFD; (*aktu&#xFFFD; (*aktu&#xFFFD; (*aktu&#xFFFD; (*aktu&#xFFFD; (*aktu&#xFFFD; (*aktu&#xFFFD; (*aktu&#xFFFD; (*aktu&#xFFFD; (*aktu&#xFFFD; (*aktu&#xFFFD; (*aktu&#xFFFD; (*aktu&#xFFFD; (*aktu&#xFFFD; (*aktu&#xFFFD; (*aktu&#xFFFD; (*aktu&#xFFFD; (*aktu&#xFFFD; (*aktu&#xFFFD; (*aktu&#xFFFD; (*aktu&#xFFFD; (*aktu&#xFFFD; (*aktu&#xFFFD; (*aktu&#xFFFD; (*aktu&#xFFFD; (*aktu&#xFFFD; (*aktu&#xFFFD; (*aktu&#xFFFD; (*aktu&#xFFFD; (*aktu&#xFFFD; (*aktu&#xFFFD; (*aktu&#xFFFD; (*aktu&#xFFFD; (*aktu&#xFFFD; (*aktu&#xFFFD; (*aktu&#xFFFD; (*aktu&#xFFFD; (*aktu&#xFFFD; (*aktu&#xFFFD; (*aktu&#xFFFD; (*aktu&#xFFFD; (*aktu&#xFFFD; (*aktu&#xFFFD; (*aktu&#xFFFD; (*aktu&#xFFFD; (*aktu&#xFFFD; (*aktu&#xFFFD; (*aktu&#xFFFD; (*aktu&#xFFFD; (*aktu&#xFFFD; (*aktu&#xFFFD; (*aktu&#xFFFD; (*aktu&#xFFFD; (*aktu&#xFFFD; (*aktu&#xFFFD; (*aktu&#xFFFD; (*aktu&#xFFFD; (*aktu&#xFFFD; (*aktu&#xFFFD; (*aktu&#xFFFD; (*aktu&#xFFFD; (*aktu&#xFFFD; (*aktu&#xFFFD; (*aktu&#xFFFD; (*aktu&#xFFFD; (*aktu&#xFFFD; (*aktu&#xFFFD; (*aktu&#xFFFD; (*aktu&#xFFFD; (*aktu&#xFFFD; (*aktu&#xFFFD; (*aktu&#xFFFD; (*aktu&#xFFFD; (*aktu&#xFFFD; (*aktu&#xFFFD; (*aktu&#xFFFD; (*aktu&#xFFFD; (*aktu&#xFFFD; (*aktu&#xFFFD; (*aktu&#xFFFD; (*aktu&#xFFFD; (*aktu&#xFFFD; (*aktu&#xFFFD; (*aktu&#xFFFD; (*aktu&#xFFFD; (*aktu&#xFFFD; (*aktu&#xFFFD; (*aktu&#xFFFD; (*aktu&#xFFFD; (*aktu&#xFFFD; (*aktu&#xFFFD; (*aktu&#xFFFD; (*aktu&#xFFFD; (*aktu&#xFFFD; (*aktu&#xFFFD; (*aktu&#xFFFD; (*aktu&#xFFFD; (*aktu&#xFFFD; (*aktu&#xFFFD; (*aktu&#xFFFD; (*aktu&#xFFFD; (*aktu&#xFFFD; (*aktu&#xFFFD; (*aktu&#xFFFD; (*aktu&#xFFFD; (*aktu&#xFFFD; (*aktu&#xFFFD; (*aktu&#xFFFD; (*aktu&#xFFFD; (*aktu&#xFFFD; (*aktu&#xFFFD; (*aktu&#xFFFD; (*aktu&#xFFFD; (*aktu&#xFFFD; (*aktu&#xFFFD; (*aktu&#xFFFD; (*aktu&#xFFFD; (*aktu&#xFFFD; (*aktu&#xFFFD; (*aktu&#xFFFD; (*aktu&#xFFFD; (*aktu&#xFFFD; (*aktu&#xFFFD; (*aktu&#xFFFD; (*aktu&#xFFFD; (*aktu&#xFFFD; (*aktu&#xFFFD; (*aktu&#xFFFD; (*aktu&#xFFFD; (*aktu&#xFFFD; (*aktu&#xFFFD; (*aktu&#xFFFD; (*aktu&#xFFFD; (*aktu&#xFFFD; (*aktu&#xFFFD; (*aktu&#xFFFD; (*aktu&#xFFFD; (*aktu&#xFFFD; (*aktu&#xFFFD; (*aktu&#xFFFD; (*aktu&#xFFFD; (*aktu&#xFFFD; (*aktu&#xFFFD; (*aktu&#xFFFD; (*aktu&#xFFFD; (*aktu&#xFFFD; (*aktu&#xFFFD; (*aktu&#xFFFD; (*aktu&#xFFFD; (*aktu&#xFFFD; (*aktu&#xFFFD; (*aktu&#xFFFD; (*aktu&#xFFFD; (*aktu&#xFFFD; (*aktu&#xFFFD; (*aktu&#xFFFD; (*aktu&#xFFFD; (*aktu&#xFFFD; (*aktu&#xFFFD; (*aktu&#xFFFD; (*aktu&#xFFFD; (*aktu&#xFFFD; (*aktu&#xFFFD; (*aktu&#xFFFD; (*aktu&#xFFFD; (*aktu&#xFFFD; (*aktu&#xFFFD; (*aktu&#xFFFD; (*aktu&#xFFFD; (*aktu&#xFFFD; (*aktu&#xFFFD; (*aktu&#xFFFD; (*aktu&#xFFFD; (*aktu&#xFFFD; (*aktu&#xFFFD; (*aktu&#xFFFD; (*aktu&#xFFFD; (*aktu&#xFFFD; (*aktu&#xFFFD; (*aktu&#xFFFD; (*aktu&#xFFFD; (*aktu&#xFFFD; (*aktu&#xFFFD; (*aktu&#xFFFD; (*aktu&#xFFFD; (*aktu&#xFFFD; (*aktu&#xFFFD; (*aktu&#xFFFD; (*aktu&#xFFFD; (*aktu&#xFFFD; (*aktu&#xFFFD; (*aktu&#xFFFD; (*aktu&#xFFFD; (*aktu&#xFFFD; (*aktu&#xFFFD; (*aktu&#xFFFD; (*aktu&#xFFFD; (*aktu&#xFFFD; (*aktu&#xFFFD; (*aktu&#xFFFD; (*aktu&#xFFFD; (*aktu&#xFFFD; (*aktu&#xFFFD; (*aktu&#xFFFD; (*aktu&#xFFFD; (*aktu&#xFFFD; (*aktu&#xFFFD; (*aktu&#xFFFD; (*aktu&#xFFFD; (*aktu&#xFFFD; (*aktu&#xFFFD; (*aktu&#xFFFD; (*aktu&#xFFFD; (*aktu&#xFFFD; (*aktu&#xFFFD; (*aktu&#xFFFD; (*aktu&#xFFFD; (*aktu&#xFFFD; (*aktu&#xFFFD; (*aktu&#xFFFD; (*aktu&#xFFFD; (*aktu&#xFFFD; (*aktu&#xFFFD; (*aktu&#xFFFD; (*aktu&#xFFFD; (*aktu&#xFFFD; (*aktu&#xFFFD; (*aktu&#xFFFD; (*aktu&#xFFFD; (*aktu&#xFFFD; (*aktu&#xFFFD; (*aktu&#xFFFD; (*aktu&#xFFFD; (*aktu&#xFFFD; (*aktu&#xFFFD; (*aktu&#xFFFD; (*aktu&#xFFFD; (*aktu&#xFFFD; (*aktu&#xFFFD; (*aktu&#xFFFD; (*aktu&#xFFFD; (*aktu&#xFFFD; (*aktu&#xFFFD; (*aktu&#xFFFD; (*aktu&#xFFFD; (*aktu&#xFFFD; (*aktu&#xFFFD; (*aktu&#xFFFD; (*aktu&#xFFFD; (*aktu&#xFFFD; (*aktu&#xFFFD; (*aktu&#xFFFD; (*aktu&#xFFFD; (*aktu&#xFFFD; (*aktu&#xFFFD; (*aktu&#xFFFD; (*aktu&#xFFFD; (*aktu&#xFFFD; (*aktu&#xFFFD; (*aktu&#xFFFD; (*aktu&#xFFFD; (*aktu&#xFFFD; (*aktu&#xFFFD; (*aktu&#xFFFD; (*aktu&#xFFFD; (*aktu&#xFFFD; (*aktu&#xFFFD; (*aktu&#xFFFD; (*aktu&#xFFFD; (*aktu&#xFFFD; (*aktu&#xFFFD; (*aktu&#xFFFD; (*aktu&#xFFFD; (*aktu&#xFFFD; (*aktu&#xFFFD; (*aktu&#xFFFD; (*aktu&#xFFFD; (*aktu&#xFFFD; (*aktu&#xFFFD; (*aktu&#xFFFD; (*aktu&#xFFFD; (*aktu&#xFFFD; (*aktu&#xFFFD; (*aktu&#xFFFD; (*aktu&#xFFFD; (*aktu&#xFFFD; (*aktu&#xFFFD; (*aktu&#xFFFD; (*aktu&#xFFFD; (*aktu&#xFFFD; (*aktu&#xFFFD; (*aktu&#xFFFD; (*aktu&#xFFFD; (*aktu&#xFFFD; (*aktu&#xFFFD; (*aktu&#xFFFD; (*aktu&#xFFFD; (*aktu&#xFFFD; (*aktu&#xFFFD; (*aktu&#xFFFD; (*aktu&#xFFFD; (*aktu&#xFFFD; (*aktu&#xFFFD; (*aktu&#xFFFD; (*aktu&#xFFFD; (*aktu&#xFFFD; (*aktu&#xFFFD; (*aktu&#xFFFD; (*aktu&#xFFFD; (*aktu&#xFFFD; (*aktu&#xFFFD; (*aktu&#xFFFD; (*aktu&#xFFFD; (*aktu&#xFFFD; (*aktu&#xFFFD; (*aktu&#xFFFD; (*aktu&#xFFFD; (*aktu&#xFFFD; (*aktu&#xFFFD; (*aktu&#xFFFD; (*aktu&#xFFFD; (*aktu&#xFFFD; (*aktu&#xFFFD; (*aktu&#xFFFD; (*aktu&#xFFFD; (*aktu&#xFFFD; (*aktu&#xFFFD; (*aktu&#xFFFD; (*aktu&#xFFFD; (*aktu&#xFFFD; (*aktu&#xFFFD; (*aktu&#xFFFD; (*aktu&#xFFFD; (*aktu&#xFFFD; (*aktu&#xFFFD; (*aktu&#xFFFD; (*aktu&#xFFFD; (*aktu&#xFFFD; (*aktu&#xFFFD; (*aktu&#xFFFD; (*aktu&#xFFFD; (*aktu&#xFFFD; (*aktu&#xFFFD; (*aktu&#xFFFD; (*aktu&#xFFFD; (*aktu&#xFFFD; (*aktu&#xFFFD; (*aktu&#xFFFD; (*aktu&#xFFFD; (*aktu&#xFFFD; (*aktu&#xFFFD; (*aktu&#xFFFD; (*aktu&#xFFFD; (*aktu&#xFFFD; (*aktu&#xFFFD; (*aktu&#xFFFD; (*aktu&#xFFFD; (*aktu&#xFFFD; (*aktu&#xFFFD; (*aktu&#xFFFD; (*aktu&#xFFFD; (*aktu&#xFFFD; (*aktu&#xFFFD; (*aktu&#xFFFD; (*aktu&#xFFFD; (*aktu&#xFFFD; (*aktu&#xFFFD; (*aktu&#xFFFD; (*aktu&#xFFFD; (*aktu&#xFFFD; (*aktu&#xFFFD; (*aktu&#xFFFD; (*aktu&#xFFFD; (*aktu&#xFFFD; (*aktu&#xFFFD; (*aktu&#xFFFD; (*aktu&#xFFFD; (*aktu&#xFFFD; (*aktu&#xFFFD; (*aktu&#xFFFD; (*aktu&#xFFFD; (*aktu&#xFFFD; (*aktu&#xFFFD; (*aktu&#xFFFD; (*aktu&#xFFFD; (*aktu&#xFFFD; (*aktu&#xFFFD; (*aktu&#xFFFD; (*aktu&#xFFFD; (*aktu&#xFFFD; (*aktu&#xFFFD; (*aktu&#xFFFD; (*aktu&#xFFFD; (*aktu&#xFFFD; (*aktu&#xFFFD; (*aktu&#xFFFD; (*aktu&#xFFFD; (*aktu&#xFFFD; (*aktu&#xFFFD; (*aktu&#xFFFD; (*aktu&#xFFFD; (*aktu&#xFFFD; (*aktu&#xFFFD; (*aktu&#xFFFD; (*aktu&#xFFFD; (*aktu&#xFFFD; (*aktu&#xFFFD; (*aktu&#xFFFD; (*aktu&#xFFFD; (*aktu&#xFFFD; (*aktu&#xFFFD; (*aktu&#xFFFD; (*aktu&#xFFFD; (*aktu&#xFFFD; (*aktu&#xFFFD; (*aktu&#xFFFD; (*aktu&#xFFFD; (*aktu&#xFFFD; (*aktu&#xFFFD; (*aktu&#xFFFD; (*aktu&#xFFFD; (*aktu&#xFFFD; (*aktu&#xFFFD; (*aktu&#xFFFD; (*aktu&#xFFFD; (*aktu&#xFFFD; (*aktu&#xFFFD; (*aktu&#xFFFD; (*aktu&#xFFFD; (*aktu&#xFFFD; (*aktu&#xFFFD; (*aktu&#xFFFD; (*aktu&#xFFFD; (*aktu&#xFFFD; (*aktu&#xFFFD; (*aktu&#xFFFD; (*aktu&#xFFFD; (*aktu&#xFFFD; (*aktu&#xFFFD; (*aktu&#xFFFD; (*aktu&#xFFFD; (*aktu&#xFFFD; (*aktu&#xFFFD; (*aktu&#xFFFD; (*aktu&#xFFFD; (*aktu&#xFFFD; (*aktu&#xFFFD; (*aktu&#xFFFD; (*aktu&#xFFFD; (*aktu&#xFFFD; (*aktu&#xFFFD; (*aktu&#xFFFD; (*aktu&#xFFFD; (*aktu&#xFFFD; (*aktu&#xFFFD; (*aktu&#xFFFD; (*aktu&#xFFFD; (*aktu&#xFFFD; (*aktu&#xFFFD; (*aktu&#xFFFD; (*aktu&#xFFFD; (*aktu&#xFFFD; (*aktu&#xFFFD; (*aktu&#xFFFD; (*aktu&#xFFFD; (*aktu&#xFFFD; (*aktu&#xFFFD; (*aktu&#xFFFD; (*aktu&#xFFFD; (*aktu&#xFFFD; (*aktu&#xFFFD; (*aktu&#xFFFD; (*aktu&#xFFFD; (*aktu&#xFFFD; (*aktu&#xFFFD; (*aktu&#xFFFD; (*aktu&#xFFFD; (*aktu&#xFFFD; (*aktu&#xFFFD; (*aktu&#xFFFD; (*aktu&#xFFFD; (*aktu&#xFFFD; (*aktu&#xFFFD; (*aktu&#xFFFD; (*aktu&#xFFFD; (*aktu&#xFFFD; (*aktu&#xFFFD; (*aktu&#xFFFD; (*aktu&#xFFFD; (*aktu&#xFFFD; (*aktu&#xFFFD; (*aktu&#xFFFD; (*aktu&#xFFFD; (*aktu&#xFFFD; (*aktu&#xFFFD; (*aktu&#xFFFD; (*aktu&#xFFFD; (*aktu&#xFFFD; (*aktu&#xFFFD; (*aktu&#xFFFD; (*aktu&#xFFFD; (*aktu&#xFFFD; (*aktu&#xFFFD; (*aktu&#xFFFD; (*aktu&#xFFFD; (*aktu&#xFFFD; (*aktu&#xFFFD; (*aktu&#xFFFD; (*aktu&#xFFFD; (*aktu&#xFFFD; (*aktu&#xFFFD; (*aktu&#xFFFD; (*aktu&#xFFFD; (*aktu&#xFFFD; (*aktu&#xFFFD; (*aktu&#xFFFD; (*aktu&#xFFFD; (*aktu&#xFFFD; (*aktu&#xFFFD; (*aktu&#xFFFD; (*aktu&#xFFFD; (*aktu&#xFFFD; (*aktu&#xFFFD; (*aktu&#xFFFD; (*aktu&#xFFFD; (*aktu&#xFFFD; (*aktu&#xFFFD; (*aktu&#xFFFD; (*aktu&#xFFFD; (*aktu&#xFFFD; (*aktu&#xFFFD; (*aktu&#xFFFD; (*aktu&#xFFFD; (*aktu&#xFFFD; (*aktu&#xFFFD; (*aktu&#xFFFD; (*aktu&#xFFFD; (*aktu&#xFFFD; (*aktu&#xFFFD; (*aktu&#xFFFD; (*aktu&#xFFFD; (*aktu&#xFFFD; (*aktu&#xFFFD; (*aktu&#xFFFD; (*aktu&#xFFFD; (*aktu&#xFFFD; (*aktu&#xFFFD; (*aktu&#xFFFD; (*aktu&#xFFFD; (*aktu&#xFFFD; (*aktu&#xFFFD; (*aktu&#xFFFD; (*aktu&#xFFFD; (*aktu&#xFFFD; (*aktu&#xFFFD; (*aktu&#xFFFD; (*aktu&#xFFFD; (*aktu&#xFFFD; (*aktu&#xFFFD; (*aktu&#xFFFD; (*aktu&#xFFFD; (*aktu&#xFFFD; (*aktu&#xFFFD; (*aktu&#xFFFD; (*aktu&#xFFFD; (*aktu&#xFFFD; (*aktu&#xFFFD; (*aktu&#xFFFD; (*aktu&#xFFFD; (*aktu&#xFFFD; (*aktu&#xFFFD; (*aktu&#xFFFD; (*aktu&#xFFFD; (*aktu&#xFFFD; (*aktu&#xFFFD; (*aktu&#xFFFD; (*aktu&#xFFFD; (*aktu&#xFFFD; (*aktu&#xFFFD; (*aktu&#xFFFD; (*aktu&#xFFFD; (*aktu&#xFFFD; (*aktu&#xFFFD; (*aktu&#xFFFD; (*aktu&#xFFFD; (*aktu&#xFFFD; (*aktu&#xFFFD; (*aktu&#xFFFD; (*aktu&#xFFFD; (*aktu&#xFFFD; (*aktu&#xFFFD; (*aktu&#xFFFD; (*aktu&#xFFFD; (*aktu&#xFFFD; (*aktu&#xFFFD; (*aktu&#xFFFD; (*aktu&#xFFFD; (*aktu&#xFFFD; (*aktu&#xFFFD; (*aktu&#xFFFD; (*aktu&#xFFFD; (*aktu&#xFFFD; (*aktu&#xFFFD; (*aktu&#xFFFD; (*aktu&#xFFFD; (*aktu&#xFFFD; (*aktu&#xFFFD; (*aktu&#xFFFD; (*aktu&#xFFFD; (*aktu&#xFFFD; (*aktu&#xFFFD; (*aktu&#xFFFD; (*aktu&#xFFFD; (*aktu&#xFFFD; (*aktu&#xFFFD; (*aktu&#xFFFD; (*aktu&#xFFFD; (*aktu&#xFFFD; (*aktu&#xFFFD; (*aktu&#xFFFD; (*aktu&#xFFFD; (*aktu&#xFFFD; (*aktu&#xFFFD; (*aktu&#xFFFD; (*aktu&#xFFFD; (*aktu&#xFFFD; (*aktu&#xFFFD; (*aktu&#xFFFD; (*aktu&#xFFFD; (*aktu&#xFFFD; (*aktu&#xFFFD; (*aktu&#xFFFD; (*aktu&#xFFFD; (*aktu&#xFFFD; (*aktu&#xFFFD; (*aktu&#xFFFD; (*aktu&#xFFFD; (*aktu&#xFFFD; (*aktu&#xFFFD; (*aktu&#xFFFD; (*aktu&#xFFFD; (*aktu&#xFFFD; (*aktu&#xFFFD; (*aktu&#xFFFD; (*aktu&#xFFFD; (*aktu&#xFFFD; (*aktu&#xFFFD; (*aktu&#xFFFD; (*aktu&#xFFFD; (*aktu&#xFFFD; (*aktu&#xFFFD; (*aktu&#xFFFD; (*aktu&#xFFFD; (*aktu&#xFFFD; (*aktu&#xFFFD; (*aktu&#xFFFD; (*aktu&#xFFFD; (*aktu&#xFFFD; (*aktu&#xFFFD; (*aktu&#xFFFD; (*aktu&#xFFFD; (*aktu&#xFFFD; (*aktu&#xFFFD; (*aktu&#xFFFD; (*aktu&#xFFFD; (*aktu&#xFFFD; (*aktu&#xFFFD; (*aktu&#xFFFD; (*aktu&#xFFFD; (*aktu&#xFFFD; (*aktu&#xFFFD; (*aktu&#xFFFD; (*aktu&#xFFFD; (*aktu&#xFFFD; (*aktu&#xFFFD; (*aktu&#xFFFD; (*aktu&#xFFFD; (*aktu&#xFFFD; (*aktu&#xFFFD; (*aktu&#xFFFD; (*aktu&#xFFFD; (*aktu&#xFFFD; (*aktu&#xFFFD; (*aktu&#xFFFD; (*aktu&#xFFFD; (*aktu&#xFFFD; (*aktu&#xFFFD; (*aktu&#xFFFD; (*aktu&#xFFFD; (*aktu&#xFFFD; (*aktu&#xFFFD; (*aktu&#xFFFD; (*aktu&#xFFFD; (*aktu&#xFFFD; (*aktu&#xFFFD; (*aktu&#xFFFD; (*aktu&#xFFFD; (*aktu&#xFFFD; (*aktu&#xFFFD; (*aktu&#xFFFD; (*aktu&#xFFFD; (*aktu&#xFFFD; (*aktu&#xFFFD; (*aktu&#xFFFD; (*aktu&#xFFFD; (*aktu&#xFFFD; (*aktu&#xFFFD; (*aktu&#xFFFD; (*aktu&#xFFFD; (*aktu&#xFFFD; (*aktu&#xFFFD; (*aktu&#xFFFD; (*aktu&#xFFFD; (*aktu&#xFFFD; (*aktu&#xFFFD; (*aktu&#xFFFD; (*aktu&#xFFFD; (*aktu&#xFFFD; (*aktu&#xFFFD; (*aktu&#xFFFD; (*aktu&#xFFFD; (*aktu&#xFFFD; (*aktu&#xFFFD; (*aktu&#xFFFD; (*aktu&#xFFFD; (*aktu&#xFFFD; (*aktu&#xFFFD; (*aktu&#xFFFD; (*aktu&#xFFFD; (*aktu&#xFFFD; (*aktu&#xFFFD; (*aktu&#xFFFD; (*aktu&#xFFFD; (*aktu&#xFFFD; (*aktu&#xFFFD; (*aktu&#xFFFD; (*aktu&#xFFFD; (*aktu&#xFFFD; (*aktu&#xFFFD; (*aktu&#xFFFD; (*aktu&#xFFFD; (*aktu&#xFFFD; (*aktu&#xFFFD; (*aktu&#xFFFD; (*aktu&#xFFFD; (*aktu&#xFFFD; (*aktu&#xFFFD; (*aktu&#xFFFD; (*aktu&#xFFFD; (*aktu&#xFFFD; (*aktu&#xFFFD; (*aktu&#xFFFD; (*aktu&#xFFFD; (*aktu&#xFFFD; (*aktu&#xFFFD; (*aktu&#xFFFD; (*aktu&#xFFFD; (*aktu&#xFFFD; (*aktu&#xFFFD; (*aktu&#xFFFD; (*aktu&#xFFFD; (*aktu&#xFFFD; (*aktu&#xFFFD; (*aktu&#xFFFD; (*aktu&#xFFFD; (*aktu&#xFFFD; (*aktu&#xFFFD; (*aktu&#xFFFD; (*aktu&#xFFFD; (*aktu&#xFFFD; (*aktu&#xFFFD; (*aktu&#xFFFD; (*aktu&#xFFFD; (*aktu&#xFFFD; (*aktu&#xFFFD; (*aktu&#xFFFD; (*aktu&#xFFFD; (*aktu&#xFFFD; (*aktu&#xFFFD; (*aktu&#xFFFD; (*aktu&#xFFFD; (*aktu&#xFFFD; (*aktu&#xFFFD; (*aktu&#xFFFD; (*aktu&#xFFFD; (*aktu&#xFFFD; (*aktu&#xFFFD; (*aktu&#xFFFD; (*aktu&#xFFFD; (*aktu&#xFFFD; (*aktu&#xFFFD; (*aktu&#xFFFD; (*aktu&#xFFFD; (*aktu&#xFFFD; (*aktu&#xFFFD; (*aktu&#xFFFD; (*aktu&#xFFFD; (*aktu&#xFFFD; (*aktu&#xFFFD; (*aktu&#xFFFD; (*aktu&#xFFFD; (*aktu&#xFFFD; (*aktu&#xFFFD; (*aktu&#xFFFD; (*aktu&#xFFFD; (*aktu&#xFFFD; (*aktu&#xFFFD; (*aktu&#xFFFD; (*aktu&#xFFFD; (*aktu&#xFFFD; (*aktu&#xFFFD; (*aktu&#xFFFD; (*aktu&#xFFFD; (*aktu&#xFFFD; (*aktu&#xFFFD; (*aktu&#xFFFD; (*aktu&#xFFFD; (*aktu&#xFFFD; (*aktu&#xFFFD; (*aktu&#xFFFD; (*aktu&#xFFFD; (*aktu&#xFFFD; (*aktu&#xFFFD; (*aktu&#xFFFD; (*aktu&#xFFFD; (*aktu&#xFFFD; (*aktu&#xFFFD; (*aktu&#xFFFD; (*aktu&#xFFFD; (*aktu&#xFFFD; (*aktu&#xFFFD; (*aktu&#xFFFD; (*aktu&#xFFFD; (*aktu&#xFFFD; (*aktu&#xFFFD; (*aktu&#xFFFD; (*aktu&#xFFFD; (*aktu&#xFFFD; (*aktu&#xFFFD; (*aktu&#xFFFD; (*aktu&#xFFFD; (*aktu&#xFFFD; (*aktu&#xFFFD; (*aktu&#xFFFD; (*aktu&#xFFFD; (*aktu&#xFFFD; (*aktu&#xFFFD; (*aktu&#xFFFD; (*aktu&#xFFFD; (*aktu&#xFFFD; (*aktu&#xFFFD; (*aktu&#xFFFD; (*aktu&#xFFFD; (*aktu&#xFFFD; (*aktu&#xFFFD; (*aktu&#xFFFD; (*aktu&#xFFFD; (*aktu&#xFFFD; (*aktu&#xFFFD; (*aktu&#xFFFD; (*aktu&#xFFFD; (*aktu&#xFFFD; (*aktu&#xFFFD; (*aktu&#xFFFD; (*aktu&#xFFFD; (*aktu&#xFFFD; (*aktu&#xFFFD; (*aktu&#xFFFD; (*aktu&#xFFFD; (*aktu&#xFFFD; (*aktu&#xFFFD; (*aktu&#xFFFD; (*aktu&#xFFFD; (*aktu&#xFFFD; (*aktu&#xFFFD; (*aktu&#xFFFD; (*aktu&#xFFFD; (*aktu&#xFFFD; (*aktu&#xFFFD; (*aktu&#xFFFD; (*aktu&#xFFFD; (*aktu&#xFFFD; (*aktu&#xFFFD; (*aktu&#xFFFD; (*aktu&#xFFFD; (*aktu&#xFFFD; (*aktu&#xFFFD; (*aktu&#xFFFD; (*aktu&#xFFFD; (*aktu&#xFFFD; (*aktu&#xFFFD; (*aktu&#xFFFD; (*aktu&#xFFFD; (*aktu&#xFFFD; (*aktu&#xFFFD; (*aktu&#xFFFD; (*aktu&#xFFFD; (*aktu&#xFFFD; (*aktu&#xFFFD; (*aktu&#xFFFD; (*aktu&#xFFFD; (*aktu&#xFFFD; (*aktu&#xFFFD; (*aktu&#xFFFD; (*aktu&#xFFFD; (*aktu&#xFFFD; (*aktu&#xFFFD; (*aktu&#xFFFD; (*aktu&#xFFFD; (*aktu&#xFFFD; (*aktu&#xFFFD; (*aktu&#xFFFD; (*aktu&#xFFFD; (*aktu&#xFFFD; (*aktu&#xFFFD; (*aktu&#xFFFD; (*aktu&#xFFFD; (*aktu&#xFFFD; (*aktu&#xFFFD; (*aktu&#xFFFD; (*aktu&#xFFFD; (*aktu&#xFFFD; (*aktu&#xFFFD; (*aktu&#xFFFD; (*aktu&#xFFFD; (*aktu&#xFFFD; (*aktu&#xFFFD; (*aktu&#xFFFD; (*aktu&#xFFFD; (*aktu&#xFFFD; (*aktu&#xFFFD; (*aktu&#xFFFD; (*aktu&#xFFFD; (*aktu&#xFFFD; (*aktu&#xFFFD; (*aktu&#xFFFD; (*aktu&#xFFFD; (*aktu&#xFFFD; (*aktu&#xFFFD; (*aktu&#xFFFD; (*aktu&#xFFFD; (*aktu&#xFFFD; (*aktu&#xFFFD; (*aktu&#xFFFD; (*aktu&#xFFFD; (*aktu&#xFFFD; (*aktu&#xFFFD; (*aktu&#xFFFD; (*aktu&#xFFFD; (*aktu&#xFFFD; (*aktu&#xFFFD; (*aktu&#xFFFD; (*aktu&#xFFFD; (*aktu&#xFFFD; (*aktu&#xFFFD; (*aktu&#xFFFD; (*aktu&#xFFFD; (*aktu&#xFFFD; (*aktu&#xFFFD; (*aktu&#xFFFD; (*aktu&#xFFFD; (*aktu&#xFFFD; (*aktu&#xFFFD; (*aktu&#xFFFD; (*aktu&#xFFFD; (*aktu&#xFFFD; (*aktu&#xFFFD; (*aktu&#xFFFD; (*aktu&#xFFFD; (*aktu&#xFFFD; (*aktu&#xFFFD; (*aktu&#xFFFD; (*aktu&#xFFFD; (*aktu&#xFFFD; (*aktu&#xFFFD; (*aktu&#xFFFD; (*aktu&#xFFFD; (*aktu&#xFFFD; (*aktu&#xFFFD; (*aktu&#xFFFD; (*aktu&#xFFFD; (*aktu&#xFFFD; (*aktu&#xFFFD; (*aktu&#xFFFD; (*aktu&#xFFFD; (*aktu&#xFFFD; (*aktu&#xFFFD; (*aktu&#xFFFD; (*aktu&#xFFFD; (*aktu&#xFFFD; (*aktu&#xFFFD; (*aktu&#xFFFD; (*aktu&#xFFFD; (*aktu&#xFFFD; (*aktu&#xFFFD; (*aktu&#xFFFD; (*aktu&#xFFFD; (*aktu&#xFFFD; (*aktu&#xFFFD; (*aktu&#xFFFD; (*aktu&#xFFFD; (*aktu&#xFFFD; (*aktu&#xFFFD; (*aktu&#xFFFD; (*aktu&#xFFFD; (*aktu&#xFFFD; (*aktu&#xFFFD; (*aktu&#xFFFD; (*aktu&#xFFFD; (*aktu&#xFFFD; (*aktu&#xFFFD; (*aktu&#xFFFD; (*aktu&#xFFFD; (*aktu&#xFFFD; (*aktu&#xFFFD; (*aktu&#xFFFD; (*aktu&#xFFFD; (*aktu&#xFFFD; (*aktu&#xFFFD; (*aktu&#xFFFD; (*aktu&#xFFFD; (*aktu&#xFFFD; (*aktu&#xFFFD; (*aktu&#xFFFD; (*aktu&#xFFFD; (*aktu&#xFFFD; (*aktu&#xFFFD; (*aktu&#xFFFD; (*aktu&#xFFFD; (*aktu&#xFFFD; (*aktu&#xFFFD; (*aktu&#xFFFD; (*aktu&#xFFFD; (*aktu&#xFFFD; (*aktu&#xFFFD; (*aktu&#xFFFD; (*aktu&#xFFFD; (*aktu&#xFFFD; (*aktu&#xFFFD; (*aktu&#xFFFD; (*aktu&#xFFFD; (*aktu&#xFFFD; (*aktu&#xFFFD; (*aktu&#xFFFD; (*aktu&#xFFFD; (*aktu&#xFFFD; (*aktu&#xFFFD; (*aktu&#xFFFD; (*aktu&#xFFFD; (*aktu&#xFFFD; (*aktu&#xFFFD; (*aktu&#xFFFD; (*aktu&#xFFFD; (*aktu&#xFFFD; (*aktu&#xFFFD; (*aktu&#xFFFD; (*aktu&#xFFFD; (*aktu&#xFFFD; (*aktu&#xFFFD; (*aktu&#xFFFD; (*aktu&#xFFFD; (*aktu&#xFFFD; (*aktu&#xFFFD; (*aktu&#xFFFD; (*aktu&#xFFFD; (*aktu&#xFFFD; (*aktu&#xFFFD; (*aktu&#xFFFD; (*aktu&#xFFFD; (*aktu&#xFFFD; (*aktu&#xFFFD; (*aktu&#xFFFD; (*aktu&#xFFFD; (*aktu&#xFFFD; (*aktu&#xFFFD; (*aktu&#xFFFD; (*aktu&#xFFFD; (*aktu&#xFFFD; (*aktu&#xFFFD; (*aktu&#xFFFD; (*aktu&#xFFFD; (*aktu&#xFFFD; (*aktu&#xFFFD; (*aktu&#xFFFD; (*aktu&#xFFFD; (*aktu&#xFFFD; (*aktu&#xFFFD; (*aktu&#xFFFD; (*aktu&#xFFFD; (*aktu&#xFFFD; (*aktu&#xFFFD; (*aktu&#xFFFD; (*aktu&#xFFFD; (*aktu&#xFFFD; (*aktu&#xFFFD; (*aktu&#xFFFD; (*aktu&#xFFFD; (*aktu&#xFFFD; (*aktu&#xFFFD; (*aktu&#xFFFD; (*aktu&#xFFFD; (*aktu&#xFFFD; (*aktu&#xFFFD; (*aktu&#xFFFD; (*aktu&#xFFFD; (*aktu&#xFFFD; (*aktu&#xFFFD; (*aktu&#xFFFD; (*aktu&#xFFFD; (*aktu&#xFFFD; (*aktu&#xFFFD; (*aktu&#xFFFD; (*aktu&#xFFFD; (*aktu&#xFFFD; (*aktu&#xFFFD; (*aktu&#xFFFD; (*aktu&#xFFFD; (*aktu&#xFFFD; (*aktu&#xFFFD; (*aktu&#xFFFD; (*aktu&#xFFFD; (*aktu&#xFFFD; (*aktu&#xFFFD; (*aktu&#xFFFD; (*aktu&#xFFFD; (*aktu&#xFFFD; (*aktu&#xFFFD; (*aktu&#xFFFD; (*aktu&#xFFFD; (*aktu&#xFFFD; (*aktu&#xFFFD; (*aktu&#xFFFD; (*aktu&#xFFFD; (*aktu&#xFFFD; (*aktu&#xFFFD; (*aktu&#xFFFD; (*aktu&#xFFFD; (*aktu&#xFFFD; (*aktu&#xFFFD; (*aktu&#xFFFD; (*aktu&#xFFFD; (*aktu&#xFFFD; (*aktu&#xFFFD; (*aktu&#xFFFD; (*aktu&#xFFFD; (*aktu&#xFFFD; (*aktu&#xFFFD; (*aktu&#xFFFD; (*aktu&#xFFFD; (*aktu&#xFFFD; (*aktu&#xFFFD; (*aktu&#xFFFD; (*aktu&#xFFFD; (*aktu&#xFFFD; (*aktu&#xFFFD; (*aktu&#xFFFD; (*aktu&#xFFFD; (*aktu&#xFFFD; (*aktu&#xFFFD; (*aktu&#xFFFD; (*aktu&#xFFFD; (*aktu&#xFFFD; (*aktu&#xFFFD; (*aktu&#xFFFD; (*aktu&#xFFFD; (*aktu&#xFFFD; (*aktu&#xFFFD; (*aktu&#xFFFD; (*aktu&#xFFFD; (*aktu&#xFFFD; (*aktu&#xFFFD; (*aktu&#xFFFD; (*aktu&#xFFFD; (*aktu&#xFFFD; (*aktu&#xFFFD; (*aktu&#xFFFD; (*aktu&#xFFFD; (*aktu&#xFFFD; (*aktu&#xFFFD; (*aktu&#xFFFD; (*aktu&#xFFFD; (*aktu&#xFFFD; (*aktu&#xFFFD; (*aktu&#xFFFD; (*aktu&#xFFFD; (*aktu&#xFFFD; (*aktu&#xFFFD; (*aktu&#xFFFD; (*aktu&#xFFFD; (*aktu&#xFFFD; (*aktu&#xFFFD; (*aktu&#xFFFD; (*aktu&#xFFFD; (*aktu&#xFFFD; (*aktu&#xFFFD; (*aktu&#xFFFD; (*aktu&#xFFFD; (*aktu&#xFFFD; (*aktu&#xFFFD; (*aktu&#xFFFD; (*aktu&#xFFFD; (*aktu&#xFFFD; (*aktu&#xFFFD; (*aktu&#xFFFD; (*aktu&#xFFFD; (*aktu&#xFFFD; (*aktu&#xFFFD; (*aktu&#xFFFD; (*aktu&#xFFFD; (*aktu&#xFFFD; (*aktu&#xFFFD; (*aktu&#xFFFD; (*aktu&#xFFFD; (*aktu&#xFFFD; (*aktu&#xFFFD; (*aktu&#xFFFD; (*aktu&#xFFFD; (*aktu&#xFFFD; (*aktu&#xFFFD; (*aktu&#xFFFD; (*aktu&#xFFFD; (*aktu&#xFFFD; (*aktu&#xFFFD; (*aktu&#xFFFD; (*aktu&#xFFFD; (*aktu&#xFFFD; (*aktu&#xFFFD; (*aktu&#xFFFD; (*aktu&#xFFFD; (*aktu&#xFFFD; (*aktu&#xFFFD; (*aktu&#xFFFD; (*aktu&#xFFFD; (*aktu&#xFFFD; (*aktu&#xFFFD; (*aktu&#xFFFD; (*aktu&#xFFFD; (*aktu&#xFFFD; (*aktu&#xFFFD; (*aktu&#xFFFD; (*aktu&#xFFFD; (*aktu&#xFFFD; (*aktu&#xFFFD; (*aktu&#xFFFD; (*aktu&#xFFFD; (*aktu&#xFFFD; (*aktu&#xFFFD; (*aktu&#xFFFD; (*aktu&#xFFFD; (*aktu&#xFFFD; (*aktu&#xFFFD; (*aktu&#xFFFD; (*aktu&#xFFFD; (*aktu&#xFFFD; (*aktu&#xFFFD; (*aktu&#xFFFD; (*aktu&#xFFFD; (*aktu&#xFFFD; (*aktu&#xFFFD; (*aktu&#xFFFD; (*aktu&#xFFFD; (*aktu&#xFFFD; (*aktu&#xFFFD; (*aktu&#xFFFD; (*aktu&#xFFFD; (*aktu&#xFFFD; (*aktu&#xFFFD; (*aktu&#xFFFD; (*aktu&#xFFFD; (*aktu&#xFFFD; (*aktu&#xFFFD; (*aktu&#xFFFD; (*aktu&#xFFFD; (*aktu&#xFFFD; (*aktu&#xFFFD; (*aktu&#xFFFD; (*aktu&#xFFFD; (*aktu&#xFFFD; (*aktu&#xFFFD; (*aktu&#xFFFD; (*aktu&#xFFFD; (*aktu&#xFFFD; (*aktu&#xFFFD; (*aktu&#xFFFD; (*aktu&#xFFFD; (*aktu&#xFFFD; (*aktu&#xFFFD; (*aktu&#xFFFD; (*aktu&#xFFFD; (*aktu&#xFFFD; (*aktu&#xFFFD; (*aktu&#xFFFD; (*aktu&#xFFFD; (*aktu&#xFFFD; (*aktu&#xFFFD; (*aktu&#xFFFD; (*aktu&#xFFFD; (*aktu&#xFFFD; (*aktu&#xFFFD; (*aktu&#xFFFD; (*aktu&#xFFFD; (*aktu&#xFFFD; (*aktu&#xFFFD; (*aktu&#xFFFD; (*aktu&#xFFFD; (*aktu&#xFFFD; (*aktu&#xFFFD; (*aktu&#xFFFD; (*aktu&#xFFFD; (*aktu&#xFFFD; (*aktu&#xFFFD; (*aktu&#xFFFD; (*aktu&#xFFFD; (*aktu&#xFFFD; (*aktu&#xFFFD; (*aktu&#xFFFD; (*aktu&#xFFFD; (*aktu&#xFFFD; (*aktu&#xFFFD; (*aktu&#xFFFD; (*aktu&#xFFFD; (*aktu&#xFFFD; (*aktu&#xFFFD; (*aktu&#xFFFD; (*aktu&#xFFFD; (*aktu&#xFFFD; (*aktu&#xFFFD; (*aktu&#xFFFD; (*aktu&#xFFFD; (*aktu&#xFFFD; (*aktu&#xFFFD; (*aktu&#xFFFD; (*aktu&#xFFFD; (*aktu&#xFFFD; (*aktu&#xFFFD; (*aktu&#xFFFD; (*aktu&#xFFFD; (*aktu&#xFFFD; (*aktu&#xFFFD; (*aktu&#xFFFD; (*aktu&#xFFFD; (*aktu&#xFFFD; (*aktu&#xFFFD; (*aktu&#xFFFD; (*aktu&#xFFFD; (*aktu&#xFFFD; (*aktu&#xFFFD; (*aktu&#xFFFD; (*aktu&#xFFFD; (*aktu&#xFFFD; (*aktu&#xFFFD; (*aktu&#xFFFD; (*aktu&#xFFFD; (*aktu&#xFFFD; (*aktu&#xFFFD; (*aktu&#xFFFD; (*aktu&#xFFFD; (*aktu&#xFFFD; (*aktu&#xFFFD; (*aktu&#xFFFD; (*aktu&#xFFFD; (*aktu&#xFFFD; (*aktu&#xFFFD; (*aktu&#xFFFD; (*aktu&#xFFFD; (*aktu&#xFFFD; (*aktu&#xFFFD; (*aktu&#xFFFD; (*aktu&#xFFFD; (*aktu&#xFFFD; (*aktu&#xFFFD; (*aktu&#xFFFD; (*aktu&#xFFFD; (*aktu&#xFFFD; (*aktu&#xFFFD; (*aktu&#xFFFD; (*aktu&#xFFFD; (*aktu&#xFFFD; (*aktu&#xFFFD; (*aktu&#xFFFD; (*aktu&#xFFFD; (*aktu&#xFFFD; (*aktu&#xFFFD; (*aktu&#xFFFD; (*aktu&#xFFFD; (*aktu&#xFFFD; (*aktu&#xFFFD; (*aktu&#xFFFD; (*aktu&#xFFFD; (*aktu&#xFFFD; (*aktu&#xFFFD; (*aktu&#xFFFD; (*aktu&#xFFFD; (*aktu&#xFFFD; (*aktu&#xFFFD; (*aktu&#xFFFD; (*aktu&#xFFFD; (*aktu&#xFFFD; (*aktu&#xFFFD; (*aktu&#xFFFD; (*aktu&#xFFFD; (*aktu&#xFFFD; (*aktu&#xFFFD; (*aktu&#xFFFD; (*aktu&#xFFFD; (*aktu&#xFFFD; (*aktu&#xFFFD; (*aktu&#xFFFD; (*aktu&#xFFFD; (*aktu&#xFFFD; (*aktu&#xFFFD; (*aktu&#xFFFD; (*aktu&#xFFFD; (*aktu&#xFFFD; (*aktu&#xFFFD; (*aktu&#xFFFD; (*aktu&#xFFFD; (*aktu&#xFFFD; (*aktu&#xFFFD; (*aktu&#xFFFD; (*aktu&#xFFFD; (*aktu&#xFFFD; (*aktu&#xFFFD; (*aktu&#xFFFD; (*aktu&#xFFFD; (*aktu&#xFFFD; (*aktu&#xFFFD; (*aktu&#xFFFD; (*aktu&#xFFFD; (*aktu&#xFFFD; (*aktu&#xFFFD; (*aktu&#xFFFD; (*aktu&#xFFFD; (*aktu&#xFFFD; (*aktu&#xFFFD; (*aktu&#xFFFD; (*aktu&#xFFFD; (*aktu&#xFFFD; (*aktu&#xFFFD; (*aktu&#xFFFD; (*aktu&#xFFFD; (*aktu&#xFFFD; (*aktu&#xFFFD; (*aktu&#xFFFD; (*aktu&#xFFFD; (*aktu&#xFFFD; (*aktu&#xFFFD; (*aktu&#xFFFD; (*aktu&#xFFFD; (*aktu&#xFFFD; (*aktu&#xFFFD; (*aktu&#xFFFD; (*aktu&#xFFFD; (*aktu&#xFFFD; (*aktu&#xFFFD; (*aktu&#xFFFD; (*aktu&#xFFFD; (*aktu&#xFFFD; (*aktu&#xFFFD; (*aktu&#xFFFD; (*aktu&#xFFFD; (*aktu&#xFFFD; (*aktu&#xFFFD; (*aktu&#xFFFD; (*aktu&#xFFFD; (*aktu&#xFFFD; (*aktu&#xFFFD; (*aktu&#xFFFD; (*aktu&#xFFFD; (*aktu&#xFFFD; (*aktu&#xFFFD; (*aktu&#xFFFD; (*aktu&#xFFFD; (*aktu&#xFFFD; (*aktu&#xFFFD; (*aktu&#xFFFD; (*aktu&#xFFFD; (*aktu&#xFFFD; (*aktu&#xFFFD; (*aktu&#xFFFD; (*aktu&#xFFFD; (*aktu&#xFFFD; (*aktu&#xFFFD; (*aktu&#xFFFD; (*aktu&#xFFFD; (*aktu&#xFFFD; (*aktu&#xFFFD; (*aktu&#xFFFD; (*aktu&#xFFFD; (*aktu&#xFFFD; (*aktu&#xFFFD; (*aktu&#xFFFD; (*aktu&#xFFFD; (*aktu&#xFFFD; (*aktu&#xFFFD; (*aktu&#xFFFD; (*aktu&#xFFFD; (*aktu&#xFFFD; (*aktu&#xFFFD; (*aktu&#xFFFD; (*aktu&#xFFFD; (*aktu&#xFFFD; (*aktu&#xFFFD; (*aktu&#xFFFD; (*aktu&#xFFFD; (*aktu&#xFFFD; (*aktu&#xFFFD; (*aktu&#xFFFD; (*aktu&#xFFFD; (*aktu&#xFFFD; (*aktu&#xFFFD; (*aktu&#xFFFD; (*aktu&#xFFFD; (*aktu&#xFFFD; (*aktu&#xFFFD; (*aktu&#xFFFD; (*aktu&#xFFFD; (*aktu&#xFFFD; (*aktu&#xFFFD; (*aktu&#xFFFD; (*aktu&#xFFFD; (*aktu&#xFFFD; (*aktu&#xFFFD; (*aktu&#xFFFD; (*aktu&#xFFFD; (*aktu&#xFFFD; (*aktu&#xFFFD; (*aktu&#xFFFD; (*aktu&#xFFFD; (*aktu&#xFFFD; (*aktu&#xFFFD; (*aktu&#xFFFD; (*aktu&#xFFFD; (*aktu&#xFFFD; (*aktu&#xFFFD; (*aktu&#xFFFD; (*aktu&#xFFFD; (*aktu&#xFFFD; (*aktu&#xFFFD; (*aktu&#xFFFD; (*aktu&#xFFFD; (*aktu&#xFFFD; (*aktu&#xFFFD; (*aktu&#xFFFD; (*aktu&#xFFFD; (*aktu&#xFFFD; (*aktu&#xFFFD; (*aktu&#xFFFD; (*aktu&#xFFFD; (*aktu&#xFFFD; (*aktu&#xFFFD; (*aktu&#xFFFD; (*aktu&#xFFFD; (*aktu&#xFFFD; (*aktu&#xFFFD; (*aktu&#xFFFD; (*aktu&#xFFFD; (*aktu&#xFFFD; (*aktu&#xFFFD; (*aktu&#xFFFD; (*aktu&#xFFFD; (*aktu&#xFFFD; (*aktu&#xFFFD; (*aktu&#xFFFD; (*aktu&#xFFFD; (*aktu&#xFFFD; (*aktu&#xFFFD; (*aktu&#xFFFD; (*aktu&#xFFFD; (*aktu&#xFFFD; (*aktu&#xFFFD; (*aktu&#xFFFD; (*aktu&#xFFFD; (*aktu&#xFFFD; (*aktu&#xFFFD; (*aktu&#xFFFD; (*aktu&#xFFFD; (*aktu&#xFFFD; (*aktu&#xFFFD; (*aktu&#xFFFD; (*aktu&#xFFFD; (*aktu&#xFFFD; (*aktu&#xFFFD; (*aktu&#xFFFD; (*aktu&#xFFFD; (*aktu&#xFFFD; (*aktu&#xFFFD; (*aktu&#xFFFD; (*aktu&#xFFFD; (*aktu&#xFFFD; (*aktu&#xFFFD; (*aktu&#xFFFD; (*aktu&#xFFFD; (*aktu&#xFFFD; (*aktu&#xFFFD; (*aktu&#xFFFD; (*aktu&#xFFFD; (*aktu&#xFFFD; (*aktu&#xFFFD; (*aktu&#xFFFD; (*aktu&#xFFFD; (*aktu&#xFFFD; (*aktu&#xFFFD; (*aktu&#xFFFD; (*aktu&#xFFFD; (*aktu&#xFFFD; (*aktu&#xFFFD; (*aktu&#xFFFD; (*aktu&#xFFFD; (*aktu&#xFFFD; (*aktu&#xFFFD; (*aktu&#xFFFD; (*aktu&#xFFFD; (*aktu&#xFFFD; (*aktu&#xFFFD; (*aktu&#xFFFD; (*aktu&#xFFFD; (*aktu&#xFFFD; (*aktu&#xFFFD; (*aktu&#xFFFD; (*aktu&#xFFFD; (*aktu&#xFFFD; (*aktu&#xFFFD; (*aktu&#xFFFD; (*aktu&#xFFFD; (*aktu&#xFFFD; (*aktu&#xFFFD; (*aktu&#xFFFD; (*aktu&#xFFFD; (*aktu&#xFFFD; (*aktu&#xFFFD; (*aktu&#xFFFD; (*aktu&#xFFFD; (*aktu&#xFFFD; (*aktu&#xFFFD; (*aktu&#xFFFD; (*aktu&#xFFFD; (*aktu&#xFFFD; (*aktu&#xFFFD; (*aktu&#xFFFD; (*aktu&#xFFFD; (*aktu&#xFFFD; (*aktu&#xFFFD; (*aktu&#xFFFD; (*aktu&#xFFFD; (*aktu&#xFFFD; (*aktu&#xFFFD; (*aktu&#xFFFD; (*aktu&#xFFFD; (*aktu&#xFFFD; (*aktu&#xFFFD; (*aktu&#xFFFD; (*aktu&#xFFFD; (*aktu&#xFFFD; (*aktu&#xFFFD; (*aktu&#xFFFD; (*aktu&#xFFFD; (*aktu&#xFFFD; (*aktu&#xFFFD; (*aktu&#xFFFD; (*aktu&#xFFFD; (*aktu&#xFFFD; (*aktu&#xFFFD; (*aktu&#xFFFD; (*aktu&#xFFFD; (*aktu&#xFFFD; (*aktu&#xFFFD; (*aktu&#xFFFD; (*aktu&#xFFFD; (*aktu&#xFFFD; (*aktu&#xFFFD; (*aktu&#xFFFD; (*aktu&#xFFFD; (*aktu&#xFFFD; (*aktu&#xFFFD; (*aktu&#xFFFD; (*aktu&#xFFFD; (*aktu&#xFFFD; (*aktu&#xFFFD; (*aktu&#xFFFD; (*aktu&#xFFFD; (*aktu&#xFFFD; (*aktu&#xFFFD; (*aktu&#xFFFD; (*aktu&#xFFFD; (*aktu&#xFFFD; (*aktu&#xFFFD; (*aktu&#xFFFD; (*aktu&#xFFFD; (*aktu&#xFFFD; (*aktu&#xFFFD; (*aktu&#xFFFD; (*aktu&#xFFFD; (*aktu&#xFFFD; (*aktu&#xFFFD; (*aktu&#xFFFD; (*aktu&#xFFFD; (*aktu&#xFFFD; (*aktu&#xFFFD; (*aktu&#xFFFD; (*aktu&#xFFFD; (*aktu&#xFFFD; (*aktu&#xFFFD; (*aktu&#xFFFD; (*aktu&#xFFFD; (*aktu&#xFFFD; (*aktu&#xFFFD; (*aktu&#xFFFD; (*aktu&#xFFFD; (*aktu&#xFFFD; (*aktu&#xFFFD; (*aktu&#xFFFD; (*aktu&#xFFFD; (*aktu&#xFFFD; (*aktu&#xFFFD; (*aktu&#xFFFD; (*aktu&#xFFFD; (*aktu&#xFFFD; (*aktu&#xFFFD; (*aktu&#xFFFD; (*aktu&#xFFFD; (*aktu&#xFFFD; (*aktu&#xFFFD; (*aktu&#xFFFD; (*aktu&#xFFFD; (*aktu&#xFFFD; (*aktu&#xFFFD; (*aktu&#xFFFD; (*aktu&#xFFFD; (*aktu&#xFFFD; (*aktu&#xFFFD; (*aktu&#xFFFD; (*aktu&#xFFFD; (*aktu&#xFFFD; (*aktu&#xFFFD; (*aktu&#xFFFD; (*aktu&#xFFFD; (*aktu&#xFFFD; (*aktu&#xFFFD; (*aktu&#xFFFD; (*aktu&#xFFFD; (*aktu&#xFFFD; (*aktu&#xFFFD; (*aktu&#xFFFD; (*aktu&#xFFFD; (*aktu&#xFFFD; (*aktu&#xFFFD; (*aktu&#xFFFD; (*aktu&#xFFFD; (*aktu&#xFFFD; (*aktu&#xFFFD; (*aktu&#xFFFD; (*aktu&#xFFFD; (*aktu&#xFFFD; (*aktu&#xFFFD; (*aktu&#xFFFD; (*aktu&#xFFFD; (*aktu&#xFFFD; (*aktu&#xFFFD; (*aktu&#xFFFD; (*aktu&#xFFFD; (*aktu&#xFFFD; (*aktu&#xFFFD; (*aktu&#xFFFD; (*aktu&#xFFFD; (*aktu&#xFFFD; (*aktu&#xFFFD; (*aktu&#xFFFD; (*aktu&#xFFFD; (*aktu&#xFFFD; (*aktu&#xFFFD; (*aktu&#xFFFD; (*aktu&#xFFFD; (*aktu&#xFFFD; (*aktu&#xFFFD; (*aktu&#xFFFD; (*aktu&#xFFFD; (*aktu&#xFFFD; (*aktu&#xFFFD; (*aktu&#xFFFD; (*aktu&#xFFFD; (*aktu&#xFFFD; (*aktu&#xFFFD; (*aktu&#xFFFD; (*aktu&#xFFFD; (*aktu&#xFFFD; (*aktu&#xFFFD; (*aktu&#xFFFD; (*aktu&#xFFFD; (*aktu&#xFFFD; (*aktu&#xFFFD; (*aktu&#xFFFD; (*aktu&#xFFFD; (*aktu&#xFFFD; (*aktu&#xFFFD; (*aktu&#xFFFD; (*aktu&#xFFFD; (*aktu&#xFFFD; (*aktu&#xFFFD; (*aktu&#xFFFD; (*aktu&#xFFFD; (*aktu&#xFFFD; (*aktu&#xFFFD; (*aktu&#xFFFD; (*aktu&#xFFFD; (*aktu&#xFFFD; (*aktu&#xFFFD; (*aktu&#xFFFD; (*aktu&#xFFFD; (*aktu&#xFFFD; (*aktu&#xFFFD; (*aktu&#xFFFD; (*aktu&#xFFFD; (*aktu&#xFFFD; (*aktu&#xFFFD; (*aktu&#xFFFD; (*aktu&#xFFFD; (*aktu&#xFFFD; (*aktu&#xFFFD; (*aktu&#xFFFD; (*aktu&#xFFFD; (*aktu&#xFFFD; (*aktu&#xFFFD; (*aktu&#xFFFD; (*aktu&#xFFFD; (*aktu&#xFFFD; (*aktu&#xFFFD; (*aktu&#xFFFD; (*aktu&#xFFFD; (*aktu&#xFFFD; (*aktu&#xFFFD; (*aktu&#xFFFD; (*aktu&#xFFFD; (*aktu&#xFFFD; (*aktu&#xFFFD; (*aktu&#xFFFD; (*aktu&#xFFFD; (*aktu&#xFFFD; (*aktu&#xFFFD; (*aktu&#xFFFD; (*aktu&#xFFFD; (*aktu&#xFFFD; (*aktu&#xFFFD; (*aktu&#xFFFD; (*aktu&#xFFFD; (*aktu&#xFFFD; (*aktu&#xFFFD; (*aktu&#xFFFD; (*aktu&#xFFFD; (*aktu&#xFFFD; (*aktu&#xFFFD; (*aktu&#xFFFD; (*aktu&#xFFFD; (*aktu&#xFFFD; (*aktu&#xFFFD; (*aktu&#xFFFD; (*aktu&#xFFFD; (*aktu&#xFFFD; (*aktu&#xFFFD; (*aktu&#xFFFD; (*aktu&#xFFFD; (*aktu&#xFFFD; (*aktu&#xFFFD; (*aktu&#xFFFD; (*aktu&#xFFFD; (*aktu&#xFFFD; (*aktu&#xFFFD; (*aktu&#xFFFD; (*aktu&#xFFFD; (*aktu&#xFFFD; (*aktu&#xFFFD; (*aktu&#xFFFD; (*aktu&#xFFFD; (*aktu&#xFFFD; (*aktu&#xFFFD; (*aktu&#xFFFD; (*aktu&#xFFFD; (*aktu&#xFFFD; (*aktu&#xFFFD; (*aktu&#xFFFD; (*aktu&#xFFFD; (*aktu&#xFFFD; (*aktu&#xFFFD; (*aktu&#xFFFD; (*aktu&#xFFFD; (*aktu&#xFFFD; (*aktu&#xFFFD; (*aktu&#xFFFD; (*aktu&#xFFFD; (*aktu&#xFFFD; (*aktu&#xFFFD; (*aktu&#xFFFD; (*aktu&#xFFFD; (*aktu&#xFFFD; (*aktu&#xFFFD; (*aktu&#xFFFD; (*aktu&#xFFFD; (*aktu&#xFFFD; (*aktu&#xFFFD; (*aktu&#xFFFD; (*aktu&#xFFFD; (*aktu&#xFFFD; (*aktu&#xFFFD; (*aktu&#xFFFD; (*aktu&#xFFFD; (*aktu&#xFFFD; (*aktu&#xFFFD; (*aktu&#xFFFD; (*aktu&#xFFFD; (*aktu&#xFFFD; (*aktu&#xFFFD; (*aktu&#xFFFD; (*aktu&#xFFFD; (*aktu&#xFFFD; (*aktu&#xFFFD; (*aktu&#xFFFD; (*aktu&#xFFFD; (*aktu&#xFFFD; (*aktu&#xFFFD; (*aktu&#xFFFD; (*aktu&#xFFFD; (*aktu&#xFFFD; (*aktu&#xFFFD; (*aktu&#xFFFD; (*aktu&#xFFFD; (*aktu&#xFFFD; (*aktu&#xFFFD; (*aktu&#xFFFD; (*aktu&#xFFFD; (*aktu&#xFFFD; (*aktu&#xFFFD; (*aktu&#xFFFD; (*aktu&#xFFFD; (*aktu&#xFFFD; (*aktu&#xFFFD; (*aktu&#xFFFD; (*aktu&#xFFFD; (*aktu&#xFFFD; (*aktu&#xFFFD; (*aktu&#xFFFD; (*aktu&#xFFFD; (*aktu&#xFFFD; (*aktu&#xFFFD; (*aktu&#xFFFD; (*aktu&#xFFFD; (*aktu&#xFFFD; (*aktu&#xFFFD; (*aktu&#xFFFD; (*aktu&#xFFFD; (*aktu&#xFFFD; (*aktu&#xFFFD; (*aktu&#xFFFD; (*aktu&#xFFFD; (*aktu&#xFFFD; (*aktu&#xFFFD; (*aktu&#xFFFD; (*aktu&#xFFFD; (*aktu&#xFFFD; (*aktu&#xFFFD; (*aktu&#xFFFD; (*aktu&#xFFFD; (*aktu&#xFFFD; (*aktu&#xFFFD; (*aktu&#xFFFD; (*aktu&#xFFFD; (*aktu&#xFFFD; (*aktu&#xFFFD; (*aktu&#xFFFD; (*aktu&#xFFFD; (*aktu&#xFFFD; (*aktu&#xFFFD; (*aktu&#xFFFD; (*aktu&#xFFFD; (*aktu&#xFFFD; (*aktu&#xFFFD; (*aktu&#xFFFD; (*aktu&#xFFFD; (*aktu&#xFFFD; (*aktu&#xFFFD; (*aktu&#xFFFD; (*aktu&#xFFFD; (*aktu&#xFFFD; (*aktu&#xFFFD; (*aktu&#xFFFD; (*aktu&#xFFFD; (*aktu&#xFFFD; (*aktu&#xFFFD; (*aktu&#xFFFD; (*aktu&#xFFFD; (*aktu&#xFFFD; (*aktu&#xFFFD; (*aktu&#xFFFD; (*aktu&#xFFFD; (*aktu&#xFFFD; (*aktu&#xFFFD; (*aktu&#xFFFD; (*aktu&#xFFFD; (*aktu&#xFFFD; (*aktu&#xFFFD; (*aktu&#xFFFD; (*aktu&#xFFFD; (*aktu&#xFFFD; (*aktu&#xFFFD; (*aktu&#xFFFD; (*aktu&#xFFFD; (*aktu&#xFFFD; (*aktu&#xFFFD; (*aktu&#xFFFD; (*aktu&#xFFFD; (*aktu&#xFFFD; (*aktu&#xFFFD; (*aktu&#xFFFD; (*aktu&#xFFFD; (*aktu&#xFFFD; (*aktu&#xFFFD; (*aktu&#xFFFD; (*aktu&#xFFFD; (*aktu&#xFFFD; (*aktu&#xFFFD; (*aktu&#xFFFD; (*aktu&#xFFFD; (*aktu&#xFFFD; (*aktu&#xFFFD; (*aktu&#xFFFD; (*aktu&#xFFFD; (*aktu&#xFFFD; (*aktu&#xFFFD; (*aktu&#xFFFD; (*aktu&#xFFFD; (*aktu&#xFFFD; (*aktu&#xFFFD; (*aktu&#xFFFD; (*aktu&#xFFFD; (*aktu&#xFFFD; (*aktu&#xFFFD; (*aktu&#xFFFD; (*aktu&#xFFFD; (*aktu&#xFFFD; (*aktu&#xFFFD; (*aktu&#xFFFD; (*aktu&#xFFFD; (*aktu&#xFFFD; (*aktu&#xFFFD; (*aktu&#xFFFD; (*aktu&#xFFFD; (*aktu&#xFFFD; (*aktu&#xFFFD; (*aktu&#xFFFD; (*aktu&#xFFFD; (*aktu&#xFFFD; (*aktu&#xFFFD; (*aktu&#xFFFD; (*aktu&#xFFFD; (*aktu&#xFFFD; (*aktu&#xFFFD; (*aktu&#xFFFD; (*aktu&#xFFFD; (*aktu&#xFFFD; (*aktu&#xFFFD; (*aktu&#xFFFD; (*aktu&#xFFFD; (*aktu&#xFFFD; (*aktu&#xFFFD; (*aktu&#xFFFD; (*aktu&#xFFFD; (*aktu&#xFFFD; (*aktu&#xFFFD; (*aktu&#xFFFD; (*aktu&#xFFFD; (*aktu&#xFFFD; (*aktu&#xFFFD; (*aktu&#xFFFD; (*aktu&#xFFFD; (*aktu&#xFFFD; (*aktu&#xFFFD; (*aktu&#xFFFD; (*aktu&#xFFFD; (*aktu&#xFFFD; (*aktu&#xFFFD; (*aktu&#xFFFD; (*aktu&#xFFFD; (*aktu&#xFFFD; (*aktu&#xFFFD; (*aktu&#xFFFD; (*aktu&#xFFFD; (*aktu&#xFFFD; (*aktu&#xFFFD; (*aktu&#xFFFD; (*aktu&#xFFFD; (*aktu&#xFFFD; (*aktu&#xFFFD; (*aktu&#xFFFD; (*aktu&#xFFFD; (*aktu&#xFFFD; (*aktu&#xFFFD; (*aktu&#xFFFD; (*aktu&#xFFFD; (*aktu&#xFFFD; (*aktu&#xFFFD; (*aktu&#xFFFD; (*aktu&#xFFFD; (*aktu&#xFFFD; (*aktu&#xFFFD; (*aktu&#xFFFD; (*aktu&#xFFFD; (*aktu&#xFFFD; (*aktu&#xFFFD; (*aktu&#xFFFD; (*aktu&#xFFFD; (*aktu&#xFFFD; (*aktu&#xFFFD; (*aktu&#xFFFD; (*aktu&#xFFFD; (*aktu&#xFFFD; (*aktu&#xFFFD; (*aktu&#xFFFD; (*aktu&#xFFFD; (*aktu&#xFFFD; (*aktu&#xFFFD; (*aktu&#xFFFD; (*aktu&#xFFFD; (*aktu&#xFFFD; (*aktu&#xFFFD; (*aktu&#xFFFD; (*aktu&#xFFFD; (*aktu&#xFFFD; (*aktu&#xFFFD; (*aktu&#xFFFD; (*aktu&#xFFFD; (*aktu&#xFFFD; (*aktu&#xFFFD; (*aktu&#xFFFD; (*aktu&#xFFFD; (*aktu&#xFFFD; (*aktu&#xFFFD; (*aktu&#xFFFD; (*aktu&#xFFFD; (*aktu&#xFFFD; (*aktu&#xFFFD; (*aktu&#xFFFD; (*aktu&#xFFFD; (*aktu&#xFFFD; (*aktu&#xFFFD; (*aktu&#xFFFD; (*aktu&#xFFFD; (*aktu&#xFFFD; (*aktu&#xFFFD; (*aktu&#xFFFD; (*aktu&#xFFFD; (*aktu&#xFFFD; (*aktu&#xFFFD; (*aktu&#xFFFD; (*aktu&#xFFFD; (*aktu&#xFFFD; (*aktu&#xFFFD; (*aktu&#xFFFD; (*aktu&#xFFFD; (*aktu&#xFFFD; (*aktu&#xFFFD; (*aktu&#xFFFD; (*aktu&#xFFFD; (*aktu&#xFFFD; (*aktu&#xFFFD; (*aktu&#xFFFD; (*aktu&#xFFFD; (*aktu&#xFFFD; (*aktu&#xFFFD; (*aktu&#xFFFD; (*aktu&#xFFFD; (*aktu&#xFFFD; (*aktu&#xFFFD; (*aktu&#xFFFD; (*aktu&#xFFFD; (*aktu&#xFFFD; (*aktu&#xFFFD; (*aktu&#xFFFD; (*aktu&#xFFFD; (*aktu&#xFFFD; (*aktu&#xFFFD; (*aktu&#xFFFD; (*aktu&#xFFFD; (*aktu&#xFFFD; (*aktu&#xFFFD; (*aktu&#xFFFD; (*aktu&#xFFFD; (*aktu&#xFFFD; (*aktu&#xFFFD; (*aktu&#xFFFD; (*aktu&#xFFFD; (*aktu&#xFFFD; (*aktu&#xFFFD; (*aktu&#xFFFD; (*aktu&#xFFFD; (*aktu&#xFFFD; (*aktu&#xFFFD; (*aktu&#xFFFD; (*aktu&#xFFFD; (*aktu&#xFFFD; (*aktu&#xFFFD; (*aktu&#xFFFD; (*aktu&#xFFFD; (*aktu&#xFFFD; (*aktu&#xFFFD; (*aktu&#xFFFD; (*aktu&#xFFFD; (*aktu&#xFFFD; (*aktu&#xFFFD; (*aktu&#xFFFD; (*aktu&#xFFFD; (*aktu&#xFFFD; (*aktu&#xFFFD; (*aktu&#xFFFD; (*aktu&#xFFFD; (*aktu&#xFFFD; (*aktu&#xFFFD; (*aktu&#xFFFD; (*aktu&#xFFFD; (*aktu&#xFFFD; (*aktu&#xFFFD; (*aktu&#xFFFD; (*aktu&#xFFFD; (*aktu&#xFFFD; (*aktu&#xFFFD; (*aktu&#xFFFD; (*aktu&#xFFFD; (*aktu&#xFFFD; (*aktu&#xFFFD; (*aktu&#xFFFD; (*aktu&#xFFFD; (*aktu&#xFFFD; (*aktu&#xFFFD; (*aktu&#xFFFD; (*aktu&#xFFFD; (*aktu&#xFFFD; (*aktu&#xFFFD; (*aktu&#xFFFD; (*aktu&#xFFFD; (*aktu&#xFFFD; (*aktu&#xFFFD; (*aktu&#xFFFD; (*aktu&#xFFFD; (*aktu&#xFFFD; (*aktu&#xFFFD; (*aktu&#xFFFD; (*aktu&#xFFFD; (*aktu&#xFFFD; (*aktu&#xFFFD; (*aktu&#xFFFD; (*aktu&#xFFFD; (*aktu&#xFFFD; (*aktu&#xFFFD; (*aktu&#xFFFD; (*aktu&#xFFFD; (*aktu&#xFFFD; (*aktu&#xFFFD; (*aktu&#xFFFD; (*aktu&#xFFFD; (*aktu&#xFFFD; (*aktu&#xFFFD; (*aktu&#xFFFD; (*aktu&#xFFFD; (*aktu&#xFFFD; (*aktu&#xFFFD; (*aktu&#xFFFD; (*aktu&#xFFFD; (*aktu&#xFFFD; (*aktu&#xFFFD; (*aktu&#xFFFD; (*aktu&#xFFFD; (*aktu&#xFFFD; (*aktu&#xFFFD; (*aktu&#xFFFD; (*aktu&#xFFFD; (*aktu&#xFFFD; (*aktu&#xFFFD; (*aktu&#xFFFD; (*aktu&#xFFFD; (*aktu&#xFFFD; (*aktu&#xFFFD; (*aktu&#xFFFD; (*aktu&#xFFFD; (*aktu&#xFFFD; (*aktu&#xFFFD; (*aktu&#xFFFD; (*aktu&#xFFFD; (*aktu&#xFFFD; (*aktu&#xFFFD; (*aktu&#xFFFD; (*aktu&#xFFFD; (*aktu&#xFFFD; (*aktu&#xFFFD; (*aktu&#xFFFD; (*aktu&#xFFFD; (*aktu&#xFFFD; (*aktu&#xFFFD; (*aktu&#xFFFD; (*aktu&#xFFFD; (*aktu&#xFFFD; (*aktu&#xFFFD; (*aktu&#xFFFD; (*aktu&#xFFFD; (*aktu&#xFFFD; (*aktu&#xFFFD; (*aktu&#xFFFD; (*aktu&#xFFFD; (*aktu&#xFFFD; (*aktu&#xFFFD; (*aktu&#xFFFD; (*aktu&#xFFFD; (*aktu&#xFFFD; (*aktu&#xFFFD; (*aktu&#xFFFD; (*aktu&#xFFFD; (*aktu&#xFFFD; (*aktu&#xFFFD; (*aktu&#xFFFD; (*aktu&#xFFFD; (*aktu&#xFFFD; (*aktu&#xFFFD; (*aktu&#xFFFD; (*aktu&#xFFFD; (*aktu&#xFFFD; (*aktu&#xFFFD; (*aktu&#xFFFD; (*aktu&#xFFFD; (*aktu&#xFFFD; (*aktu&#xFFFD; (*aktu&#xFFFD; (*aktu&#xFFFD; (*aktu&#xFFFD; (*aktu&#xFFFD; (*aktu&#xFFFD; (*aktu&#xFFFD; (*aktu&#xFFFD; (*aktu&#xFFFD; (*aktu&#xFFFD; (*aktu&#xFFFD; (*aktu&#xFFFD; (*aktu&#xFFFD; (*aktu&#xFFFD; (*aktu&#xFFFD; (*aktu&#xFFFD; (*aktu&#xFFFD; (*aktu&#xFFFD; (*aktu&#xFFFD; (*aktu&#xFFFD; (*aktu&#xFFFD; (*aktu&#xFFFD; (*aktu&#xFFFD; (*aktu&#xFFFD; (*aktu&#xFFFD; (*aktu&#xFFFD; (*aktu&#xFFFD; (*aktu&#xFFFD; (*aktu&#xFFFD; (*aktu&#xFFFD; (*aktu&#xFFFD; (*aktu&#xFFFD; (*aktu&#xFFFD; (*aktu&#xFFFD; (*aktu&#xFFFD; (*aktu&#xFFFD; (*aktu&#xFFFD; (*aktu&#xFFFD; (*aktu&#xFFFD; (*aktu&#xFFFD; (*aktu&#xFFFD; (*aktu&#xFFFD; (*aktu&#xFFFD; (*aktu&#xFFFD; (*aktu&#xFFFD; (*aktu&#xFFFD; (*aktu&#xFFFD; (*aktu&#xFFFD; (*aktu&#xFFFD; (*aktu&#xFFFD; (*aktu&#xFFFD; (*aktu&#xFFFD; (*aktu&#xFFFD; (*aktu&#xFFFD; (*aktu&#xFFFD; (*aktu&#xFFFD; (*aktu&#xFFFD; (*aktu&#xFFFD; (*aktu&#xFFFD; (*aktu&#xFFFD; (*aktu&#xFFFD; (*aktu&#xFFFD; (*aktu&#xFFFD; (*aktu&#xFFFD; (*aktu&#xFFFD; (*aktu&#xFFFD; (*aktu&#xFFFD; (*aktu&#xFFFD; (*aktu&#xFFFD; (*aktu&#xFFFD; (*aktu&#xFFFD; (*aktu&#xFFFD; (*aktu&#xFFFD; (*aktu&#xFFFD; (*aktu&#xFFFD; (*aktu&#xFFFD; (*aktu&#xFFFD; (*aktu&#xFFFD; (*aktu&#xFFFD; (*aktu&#xFFFD; (*aktu&#xFFFD; (*aktu&#xFFFD; (*aktu&#xFFFD; (*aktu&#xFFFD; (*aktu&#xFFFD; (*aktu&#xFFFD; (*aktu&#xFFFD; (*aktu&#xFFFD; (*aktu&#xFFFD; (*aktu&#xFFFD; (*aktu&#xFFFD; (*aktu&#xFFFD; (*aktu&#xFFFD; (*aktu&#xFFFD; (*aktu&#xFFFD; (*aktu&#xFFFD; (*aktu&#xFFFD; (*aktu&#xFFFD; (*aktu&#xFFFD; (*aktu&#xFFFD; (*aktu&#xFFFD; (*aktu&#xFFFD; (*aktu&#xFFFD; (*aktu&#xFFFD; (*aktu&#xFFFD; (*aktu&#xFFFD; (*aktu&#xFFFD; (*aktu&#xFFFD; (*aktu&#xFFFD; (*aktu&#xFFFD; (*aktu&#xFFFD; (*aktu&#xFFFD; (*aktu&#xFFFD; (*aktu&#xFFFD; (*aktu&#xFFFD; (*aktu&#xFFFD; (*aktu&#xFFFD; (*aktu&#xFFFD; (*aktu&#xFFFD; (*aktu&#xFFFD; (*aktu&#xFFFD; (*aktu&#xFFFD; (*aktu&#xFFFD; (*aktu&#xFFFD; (*aktu&#xFFFD; (*aktu&#xFFFD; (*aktu&#xFFFD; (*aktu&#xFFFD; (*aktu&#xFFFD; (*aktu&#xFFFD; (*aktu&#xFFFD; (*aktu&#xFFFD; (*aktu&#xFFFD; (*aktu&#xFFFD; (*aktu&#xFFFD; (*aktu&#xFFFD; (*aktu&#xFFFD; (*aktu&#xFFFD; (*aktu&#xFFFD; (*aktu&#xFFFD; (*aktu&#xFFFD; (*aktu&#xFFFD; (*aktu&#xFFFD; (*aktu&#xFFFD; (*aktu&#xFFFD; (*aktu&#xFFFD; (*aktu&#xFFFD; (*aktu&#xFFFD; (*aktu&#xFFFD; (*aktu&#xFFFD; (*aktu&#xFFFD; (*aktu&#xFFFD; (*aktu&#xFFFD; (*aktu&#xFFFD; (*aktu&#xFFFD; (*aktu&#xFFFD; (*aktu&#xFFFD; (*aktu&#xFFFD; (*aktu&#xFFFD; (*aktu&#xFFFD; (*aktu&#xFFFD; (*aktu&#xFFFD; (*aktu&#xFFFD; (*aktu&#xFFFD; (*aktu&#xFFFD; (*aktu&#xFFFD; (*aktu&#xFFFD; (*aktu&#xFFFD; (*aktu&#xFFFD; (*aktu&#xFFFD; (*aktu&#xFFFD; (*aktu&#xFFFD; (*aktu&#xFFFD; (*aktu&#xFFFD; (*aktu&#xFFFD; (*aktu&#xFFFD; (*aktu&#xFFFD; (*aktu&#xFFFD; (*aktu&#xFFFD; (*aktu&#xFFFD; (*aktu&#xFFFD; (*aktu&#xFFFD; (*aktu&#xFFFD; (*aktu&#xFFFD; (*aktu&#xFFFD; (*aktu&#xFFFD; (*aktu&#xFFFD; (*aktu&#xFFFD; (*aktu&#xFFFD; (*aktu&#xFFFD; (*aktu&#xFFFD; (*aktu&#xFFFD; (*aktu&#xFFFD; (*aktu&#xFFFD; (*aktu&#xFFFD; (*aktu&#xFFFD; (*aktu&#xFFFD; (*aktu&#xFFFD; (*aktu&#xFFFD; (*aktu&#xFFFD; (*aktu&#xFFFD; (*aktu&#xFFFD; (*aktu&#xFFFD; (*aktu&#xFFFD; (*aktu&#xFFFD; (*aktu&#xFFFD; (*aktu&#xFFFD; (*aktu&#xFFFD; (*aktu&#xFFFD; (*aktu&#xFFFD; (*aktu&#xFFFD; (*aktu&#xFFFD; (*aktu&#xFFFD; (*aktu&#xFFFD; (*aktu&#xFFFD; (*aktu&#xFFFD; (*aktu&#xFFFD; (*aktu&#xFFFD; (*aktu&#xFFFD; (*aktu&#xFFFD; (*aktu&#xFFFD; (*aktu&#xFFFD; (*aktu&#xFFFD; (*aktu&#xFFFD; (*aktu&#xFFFD; (*aktu&#xFFFD; (*aktu&#xFFFD; (*aktu&#xFFFD; (*aktu&#xFFFD; (*aktu&#xFFFD; (*aktu&#xFFFD; (*aktu&#xFFFD; (*aktu&#xFFFD; (*aktu&#xFFFD; (*aktu&#xFFFD; (*aktu&#xFFFD; (*aktu&#xFFFD; (*aktu&#xFFFD; (*aktu&#xFFFD; (*aktu&#xFFFD; (*aktu&#xFFFD; (*aktu&#xFFFD; (*aktu&#xFFFD; (*aktu&#xFFFD; (*aktu&#xFFFD; (*aktu&#xFFFD; (*aktu&#xFFFD; (*aktu&#xFFFD; (*aktu&#xFFFD; (*aktu&#xFFFD; (*aktu&#xFFFD; (*aktu&#xFFFD; (*aktu&#xFFFD; (*aktu&#xFFFD; (*aktu&#xFFFD; (*aktu&#xFFFD; (*aktu&#xFFFD; (*aktu&#xFFFD; (*aktu&#xFFFD; (*aktu&#xFFFD; (*aktu&#xFFFD; (*aktu&#xFFFD; (*aktu&#xFFFD; (*aktu&#xFFFD; (*aktu&#xFFFD; (*aktu&#xFFFD; (*aktu&#xFFFD; (*aktu&#xFFFD; (*aktu&#xFFFD; (*aktu&#xFFFD; (*aktu&#xFFFD; (*aktu&#xFFFD; (*aktu&#xFFFD; (*aktu&#xFFFD; (*aktu&#xFFFD; (*aktu&#xFFFD; (*aktu&#xFFFD; (*aktu&#xFFFD; (*aktu&#xFFFD; (*aktu&#xFFFD; (*aktu&#xFFFD; (*aktu&#xFFFD; (*aktu&#xFFFD; (*aktu&#xFFFD; (*aktu&#xFFFD; (*aktu&#xFFFD; (*aktu&#xFFFD; (*aktu&#xFFFD; (*aktu&#xFFFD; (*aktu&#xFFFD; (*aktu&#xFFFD; (*aktu&#xFFFD; (*aktu&#xFFFD; (*aktu&#xFFFD; (*aktu&#xFFFD; (*aktu&#xFFFD; (*aktu&#xFFFD; (*aktu&#xFFFD; (*aktu&#xFFFD; (*aktu&#xFFFD; (*aktu&#xFFFD; (*aktu&#xFFFD; (*aktu&#xFFFD; (*aktu&#xFFFD; (*aktu&#xFFFD; (*aktu&#xFFFD; (*aktu&#xFFFD; (*aktu&#xFFFD; (*aktu&#xFFFD; (*aktu&#xFFFD; (*aktu&#xFFFD; (*aktu&#xFFFD; (*aktu&#xFFFD; (*aktu&#xFFFD; (*aktu&#xFFFD; (*aktu&#xFFFD; (*aktu&#xFFFD; (*aktu&#xFFFD; (*aktu&#xFFFD; (*aktu&#xFFFD; (*aktu&#xFFFD; (*aktu&#xFFFD; (*aktu&#xFFFD; (*aktu&#xFFFD; (*aktu&#xFFFD; (*aktu&#xFFFD; (*aktu&#xFFFD; (*aktu&#xFFFD; (*aktu&#xFFFD; (*aktu&#xFFFD; (*aktu&#xFFFD; (*aktu&#xFFFD; (*aktu&#xFFFD; (*aktu&#xFFFD; (*aktu&#xFFFD; (*aktu&#xFFFD; (*aktu&#xFFFD; (*aktu&#xFFFD; (*aktu&#xFFFD; (*aktu&#xFFFD; (*aktu&#xFFFD; (*aktu&#xFFFD; (*aktu&#xFFFD; (*aktu&#xFFFD; (*aktu&#xFFFD; (*aktu&#xFFFD; (*aktu&#xFFFD; (*aktu&#xFFFD; (*aktu&#xFFFD; (*aktu&#xFFFD; (*aktu&#xFFFD; (*aktu&#xFFFD; (*aktu&#xFFFD; (*aktu&#xFFFD; (*aktu&#xFFFD; (*aktu&#xFFFD; (*aktu&#xFFFD; (*aktu&#xFFFD; (*aktu&#xFFFD; (*aktu&#xFFFD; (*aktu&#xFFFD; (*aktu&#xFFFD; (*aktu&#xFFFD; (*aktu&#xFFFD; (*aktu&#xFFFD; (*aktu&#xFFFD; (*aktu&#xFFFD; (*aktu&#xFFFD; (*aktu&#xFFFD; (*aktu&#xFFFD; (*aktu&#xFFFD; (*aktu&#xFFFD; (*aktu&#xFFFD; (*aktu&#xFFFD; (*aktu&#xFFFD; (*aktu&#xFFFD; (*aktu&#xFFFD; (*aktu&#xFFFD; (*aktu&#xFFFD; (*aktu&#xFFFD; (*aktu&#xFFFD; (*aktu&#xFFFD; (*aktu&#xFFFD; (*aktu&#xFFFD; (*aktu&#xFFFD; (*aktu&#xFFFD; (*aktu&#xFFFD; (*aktu&#xFFFD; (*aktu&#xFFFD; (*aktu&#xFFFD; (*aktu&#xFFFD; (*aktu&#xFFFD; (*aktu&#xFFFD; (*aktu&#xFFFD; (*aktu&#xFFFD; (*aktu&#xFFFD; (*aktu&#xFFFD; (*aktu&#xFFFD; (*aktu&#xFFFD; (*aktu&#xFFFD; (*aktu&#xFFFD; (*aktu&#xFFFD; (*aktu&#xFFFD; (*aktu&#xFFFD; (*aktu&#xFFFD; (*aktu&#xFFFD; (*aktu&#xFFFD; (*aktu&#xFFFD; (*aktu&#xFFFD; (*aktu&#xFFFD; (*aktu&#xFFFD; (*aktu&#xFFFD; (*aktu&#xFFFD; (*aktu&#xFFFD; (*aktu&#xFFFD; (*aktu&#xFFFD; (*aktu&#xFFFD; (*aktu&#xFFFD; (*aktu&#xFFFD; (*aktu&#xFFFD; (*aktu&#xFFFD; (*aktu&#xFFFD; (*aktu&#xFFFD; (*aktu&#xFFFD; (*aktu&#xFFFD; (*aktu&#xFFFD; (*aktu&#xFFFD; (*aktu&#xFFFD; (*aktu&#xFFFD; (*aktu&#xFFFD; (*aktu&#xFFFD; (*aktu&#xFFFD; (*aktu&#xFFFD; (*aktu&#xFFFD; (*aktu&#xFFFD; (*aktu&#xFFFD; (*aktu&#xFFFD; (*aktu&#xFFFD; (*aktu&#xFFFD; (*aktu&#xFFFD; (*aktu&#xFFFD; (*aktu&#xFFFD; (*aktu&#xFFFD; (*aktu&#xFFFD; (*aktu&#xFFFD; (*aktu&#xFFFD; (*aktu&#xFFFD; (*aktu&#xFFFD; (*aktu&#xFFFD; (*aktu&#xFFFD; (*aktu&#xFFFD; (*aktu&#xFFFD; (*aktu&#xFFFD; (*aktu&#xFFFD; (*aktu&#xFFFD; (*aktu&#xFFFD; (*aktu&#xFFFD; (*aktu&#xFFFD; (*aktu&#xFFFD; (*aktu&#xFFFD; (*aktu&#xFFFD; (*aktu&#xFFFD; (*aktu&#xFFFD; (*aktu&#xFFFD; (*aktu&#xFFFD; (*aktu&#xFFFD; (*aktu&#xFFFD; (*aktu&#xFFFD; (*aktu&#xFFFD; (*aktu&#xFFFD; (*aktu&#xFFFD; (*aktu&#xFFFD; (*aktu&#xFFFD; (*aktu&#xFFFD; (*aktu&#xFFFD; (*aktu&#xFFFD; (*aktu&#xFFFD; (*aktu&#xFFFD; (*aktu&#xFFFD; (*aktu&#xFFFD; (*aktu&#xFFFD; (*aktu&#xFFFD; (*aktu&#xFFFD; (*aktu&#xFFFD; (*aktu&#xFFFD; (*aktu&#xFFFD; (*aktu&#xFFFD; (*aktu&#xFFFD; (*aktu&#xFFFD; (*aktu&#xFFFD; (*aktu&#xFFFD; (*aktu&#xFFFD; (*aktu&#xFFFD; (*aktu&#xFFFD; (*aktu&#xFFFD; (*aktu&#xFFFD; (*aktu&#xFFFD; (*aktu&#xFFFD; (*aktu&#xFFFD; (*aktu&#xFFFD; (*aktu&#xFFFD; (*aktu&#xFFFD; (*aktu&#xFFFD; (*aktu&#xFFFD; (*aktu&#xFFFD; (*aktu&#xFFFD; (*aktu&#xFFFD; (*aktu&#xFFFD; (*aktu&#xFFFD; (*aktu&#xFFFD; (*aktu&#xFFFD; (*aktu&#xFFFD; (*aktu&#xFFFD; (*aktu&#xFFFD; (*aktu&#xFFFD; (*aktu&#xFFFD; (*aktu&#xFFFD; (*aktu&#xFFFD; (*aktu&#xFFFD; (*aktu&#xFFFD; (*aktu&#xFFFD; (*aktu&#xFFFD; (*aktu&#xFFFD; (*aktu&#xFFFD; (*aktu&#xFFFD; (*aktu&#xFFFD; (*aktu&#xFFFD; (*aktu&#xFFFD; (*aktu&#xFFFD; (*aktu&#xFFFD; (*aktu&#xFFFD; (*aktu&#xFFFD; (*aktu&#xFFFD; (*aktu&#xFFFD; (*aktu&#xFFFD; (*aktu&#xFFFD; (*aktu&#xFFFD; (*aktu&#xFFFD; (*aktu&#xFFFD; (*aktu&#xFFFD; (*aktu&#xFFFD; (*aktu&#xFFFD; (*aktu&#xFFFD; (*aktu&#xFFFD; (*aktu&#xFFFD; (*aktu&#xFFFD; (*aktu&#xFFFD; (*aktu&#xFFFD; (*aktu&#xFFFD; (*aktu&#xFFFD; (*aktu&#xFFFD; (*aktu&#xFFFD; (*aktu&#xFFFD; (*aktu&#xFFFD; (*aktu&#xFFFD; (*aktu&#xFFFD; (*aktu&#xFFFD; (*aktu&#xFFFD; (*aktu&#xFFFD; (*aktu&#xFFFD; (*aktu&#xFFFD; (*aktu&#xFFFD; (*aktu&#xFFFD; (*aktu&#xFFFD; (*aktu&#xFFFD; (*aktu&#xFFFD; (*aktu&#xFFFD; (*aktu&#xFFFD; (*aktu&#xFFFD; (*aktu&#xFFFD; (*aktu&#xFFFD; (*aktu&#xFFFD; (*aktu&#xFFFD; (*aktu&#xFFFD; (*aktu&#xFFFD; (*aktu&#xFFFD; (*aktu&#xFFFD; (*aktu&#xFFFD; (*aktu&#xFFFD; (*aktu&#xFFFD; (*aktu&#xFFFD; (*aktu&#xFFFD; (*aktu&#xFFFD; (*aktu&#xFFFD; (*aktu&#xFFFD; (*aktu&#xFFFD; (*aktu&#xFFFD; (*aktu&#xFFFD; (*aktu&#xFFFD; (*aktu&#xFFFD; (*aktu&#xFFFD; (*aktu&#xFFFD; (*aktu&#xFFFD; (*aktu&#xFFFD; (*aktu&#xFFFD; (*aktu&#xFFFD; (*aktu&#xFFFD; (*aktu&#xFFFD; (*aktu&#xFFFD; (*aktu&#xFFFD; (*aktu&#xFFFD; (*aktu&#xFFFD; (*aktu&#xFFFD; (*aktu&#xFFFD; (*aktu&#xFFFD; (*aktu&#xFFFD; (*aktu&#xFFFD; (*aktu&#xFFFD; (*aktu&#xFFFD; (*aktu&#xFFFD; (*aktu&#xFFFD; (*aktu&#xFFFD; (*aktu&#xFFFD; (*aktu&#xFFFD; (*aktu&#xFFFD; (*aktu&#xFFFD; (*aktu&#xFFFD; (*aktu&#xFFFD; (*aktu&#xFFFD; (*aktu&#xFFFD; (*aktu&#xFFFD; (*aktu&#xFFFD; (*aktu&#xFFFD; (*aktu&#xFFFD; (*aktu&#xFFFD; (*aktu&#xFFFD; (*aktu&#xFFFD; (*aktu&#xFFFD; (*aktu&#xFFFD; (*aktu&#xFFFD; (*aktu&#xFFFD; (*aktu&#xFFFD; (*aktu&#xFFFD; (*aktu&#xFFFD; (*aktu&#xFFFD; (*aktu&#xFFFD; (*aktu&#xFFFD; (*aktu&#xFFFD; (*aktu&#xFFFD; (*aktu&#xFFFD; (*aktu&#xFFFD; (*aktu&#xFFFD; (*aktu&#xFFFD; (*aktu&#xFFFD; (*aktu&#xFFFD; (*aktu&#xFFFD; (*aktu&#xFFFD; (*aktu&#xFFFD; (*aktu&#xFFFD; (*aktu&#xFFFD; (*aktu&#xFFFD; (*aktu&#xFFFD; (*aktu&#xFFFD; (*aktu&#xFFFD; (*aktu&#xFFFD; (*aktu&#xFFFD; (*aktu&#xFFFD; (*aktu&#xFFFD; (*aktu&#xFFFD; (*aktu&#xFFFD; (*aktu&#xFFFD; (*aktu&#xFFFD; (*aktu&#xFFFD; (*aktu&#xFFFD; (*aktu&#xFFFD; (*aktu&#xFFFD; (*aktu&#xFFFD; (*aktu&#xFFFD; (*aktu&#xFFFD; (*aktu&#xFFFD; (*aktu&#xFFFD; (*aktu&#xFFFD; (*aktu&#xFFFD; (*aktu&#xFFFD; (*aktu&#xFFFD; (*aktu&#xFFFD; (*aktu&#xFFFD; (*aktu&#xFFFD; (*aktu&#xFFFD; (*aktu&#xFFFD; (*aktu&#xFFFD; (*aktu&#xFFFD; (*aktu&#xFFFD; (*aktu&#xFFFD; (*aktu&#xFFFD; (*aktu&#xFFFD; (*aktu&#xFFFD; (*aktu&#xFFFD; (*aktu&#xFFFD; (*aktu&#xFFFD; (*aktu&#xFFFD; (*aktu&#xFFFD; (*aktu&#xFFFD; (*aktu&#xFFFD; (*aktu&#xFFFD; (*aktu&#xFFFD; (*aktu&#xFFFD; (*aktu&#xFFFD; (*aktu&#xFFFD; (*aktu&#xFFFD; (*aktu&#xFFFD; (*aktu&#xFFFD; (*aktu&#xFFFD; (*aktu&#xFFFD; (*aktu&#xFFFD; (*aktu&#xFFFD; (*aktu&#xFFFD; (*aktu&#xFFFD; (*aktu&#xFFFD; (*aktu&#xFFFD; (*aktu&#xFFFD; (*aktu&#xFFFD; (*aktu&#xFFFD; (*aktu&#xFFFD; (*aktu&#xFFFD; (*aktu&#xFFFD; (*aktu&#xFFFD; (*aktu&#xFFFD; (*aktu&#xFFFD; (*aktu&#xFFFD; (*aktu&#xFFFD; (*aktu&#xFFFD; (*aktu&#xFFFD; (*aktu&#xFFFD; (*aktu&#xFFFD; (*aktu&#xFFFD; (*aktu&#xFFFD; (*aktu&#xFFFD; (*aktu&#xFFFD; (*aktu&#xFFFD; (*aktu&#xFFFD; (*aktu&#xFFFD; (*aktu&#xFFFD; (*aktu&#xFFFD; (*aktu&#xFFFD; (*aktu&#xFFFD; (*aktu&#xFFFD; (*aktu&#xFFFD; (*aktu&#xFFFD; (*aktu&#xFFFD; (*aktu&#xFFFD; (*aktu&#xFFFD; (*aktu&#xFFFD; (*aktu&#xFFFD; (*aktu&#xFFFD; (*aktu&#xFFFD; (*aktu&#xFFFD; (*aktu&#xFFFD; (*aktu&#xFFFD; (*aktu&#xFFFD; (*aktu&#xFFFD; (*aktu&#xFFFD; (*aktu&#xFFFD; (*aktu&#xFFFD; (*aktu&#xFFFD; (*aktu&#xFFFD; (*aktu&#xFFFD; (*aktu&#xFFFD; (*aktu&#xFFFD; (*aktu&#xFFFD; (*aktu&#xFFFD; (*aktu&#xFFFD; (*aktu&#xFFFD; (*aktu&#xFFFD; (*aktu&#xFFFD; (*aktu&#xFFFD; (*aktu&#xFFFD; (*aktu&#xFFFD; (*aktu&#xFFFD; (*aktu&#xFFFD; (*aktu&#xFFFD; (*aktu&#xFFFD; (*aktu&#xFFFD; (*aktu&#xFFFD; (*aktu&#xFFFD; (*aktu&#xFFFD; (*aktu&#xFFFD; (*aktu&#xFFFD; (*aktu&#xFFFD; (*aktu&#xFFFD; (*aktu&#xFFFD; (*aktu&#xFFFD; (*aktu&#xFFFD; (*aktu&#xFFFD; (*aktu&#xFFFD; (*aktu&#xFFFD; (*aktu&#xFFFD; (*aktu&#xFFFD; (*aktu&#xFFFD; (*aktu&#xFFFD; (*aktu&#xFFFD; (*aktu&#xFFFD; (*aktu&#xFFFD; (*aktu&#xFFFD; (*aktu&#xFFFD; (*aktu&#xFFFD; (*aktu&#xFFFD; (*aktu&#xFFFD; (*aktu&#xFFFD; (*aktu&#xFFFD; (*aktu&#xFFFD; (*aktu&#xFFFD; (*aktu&#xFFFD; (*aktu&#xFFFD; (*aktu&#xFFFD; (*aktu&#xFFFD; (*aktu&#xFFFD; (*aktu&#xFFFD; (*aktu&#xFFFD; (*aktu&#xFFFD; (*aktu&#xFFFD; (*aktu&#xFFFD; (*aktu&#xFFFD; (*aktu&#xFFFD; (*aktu&#xFFFD; (*aktu&#xFFFD; (*aktu&#xFFFD; (*aktu&#xFFFD; (*aktu&#xFFFD; (*aktu&#xFFFD; (*aktu&#xFFFD; (*aktu&#xFFFD; (*aktu&#xFFFD; (*aktu&#xFFFD; (*aktu&#xFFFD; (*aktu&#xFFFD; (*aktu&#xFFFD; (*aktu&#xFFFD; (*aktu&#xFFFD; (*aktu&#xFFFD; (*aktu&#xFFFD; (*aktu&#xFFFD; (*aktu&#xFFFD; (*aktu&#xFFFD; (*aktu&#xFFFD; (*aktu&#xFFFD; (*aktu&#xFFFD; (*aktu&#xFFFD; (*aktu&#xFFFD; (*aktu&#xFFFD; (*aktu&#xFFFD; (*aktu&#xFFFD; (*aktu&#xFFFD; (*aktu&#xFFFD; (*aktu&#xFFFD; (*aktu&#xFFFD; (*aktu&#xFFFD; (*aktu&#xFFFD; (*aktu&#xFFFD; (*aktu&#xFFFD; (*aktu&#xFFFD; (*aktu&#xFFFD; (*aktu&#xFFFD; (*aktu&#xFFFD; (*aktu&#xFFFD; (*aktu&#xFFFD; (*aktu&#xFFFD; (*aktu&#xFFFD; (*aktu&#xFFFD; (*aktu&#xFFFD; (*aktu&#xFFFD; (*aktu&#xFFFD; (*aktu&#xFFFD; (*aktu&#xFFFD; (*aktu&#xFFFD; (*aktu&#xFFFD; (*aktu&#xFFFD; (*aktu&#xFFFD; (*aktu&#xFFFD; (*aktu&#xFFFD; (*aktu&#xFFFD; (*aktu&#xFFFD; (*aktu&#xFFFD; (*aktu&#xFFFD; (*aktu&#xFFFD; (*aktu&#xFFFD; (*aktu&#xFFFD; (*aktu&#xFFFD; (*aktu&#xFFFD; (*aktu&#xFFFD; (*aktu&#xFFFD; (*aktu&#xFFFD; (*aktu&#xFFFD; (*aktu&#xFFFD; (*aktu&#xFFFD; (*aktu&#xFFFD; (*aktu&#xFFFD; (*aktu&#xFFFD; (*aktu&#xFFFD; (*aktu&#xFFFD; (*aktu&#xFFFD; (*aktu&#xFFFD; (*aktu&#xFFFD; (*aktu&#xFFFD; (*aktu&#xFFFD; (*aktu&#xFFFD; (*aktu&#xFFFD; (*aktu&#xFFFD; (*aktu&#xFFFD; (*aktu&#xFFFD; (*aktu&#xFFFD; (*aktu&#xFFFD; (*aktu&#xFFFD; (*aktu&#xFFFD; (*aktu&#xFFFD; (*aktu&#xFFFD; (*aktu&#xFFFD; (*aktu&#xFFFD; (*aktu&#xFFFD; (*aktu&#xFFFD; (*aktu&#xFFFD; (*aktu&#xFFFD; (*aktu&#xFFFD; (*aktu&#xFFFD; (*aktu&#xFFFD; (*aktu&#xFFFD; (*aktu&#xFFFD; (*aktu&#xFFFD; (*aktu&#xFFFD; (*aktu&#xFFFD; (*aktu&#xFFFD; (*aktu&#xFFFD; (*aktu&#xFFFD; (*aktu&#xFFFD; (*aktu&#xFFFD; (*aktu&#xFFFD; (*aktu&#xFFFD; (*aktu&#xFFFD; (*aktu&#xFFFD; (*aktu&#xFFFD; (*aktu&#xFFFD; (*aktu&#xFFFD; (*aktu&#xFFFD; (*aktu&#xFFFD; (*aktu&#xFFFD; (*aktu&#xFFFD; (*aktu&#xFFFD; (*aktu&#xFFFD; (*aktu&#xFFFD; (*aktu&#xFFFD; (*aktu&#xFFFD; (*aktu&#xFFFD; (*aktu&#xFFFD; (*aktu&#xFFFD; (*aktu&#xFFFD; (*aktu&#xFFFD; (*aktu&#xFFFD; (*aktu&#xFFFD; (*aktu&#xFFFD; (*aktu&#xFFFD; (*aktu&#xFFFD; (*aktu&#xFFFD; (*aktu&#xFFFD; (*aktu&#xFFFD; (*aktu&#xFFFD; (*aktu&#xFFFD; (*aktu&#xFFFD; (*aktu&#xFFFD; (*aktu&#xFFFD; (*aktu&#xFFFD; (*aktu&#xFFFD; (*aktu&#xFFFD; (*aktu&#xFFFD; (*aktu&#xFFFD; (*aktu&#xFFFD; (*aktu&#xFFFD; (*aktu&#xFFFD; (*aktu&#xFFFD; (*aktu&#xFFFD; (*aktu&#xFFFD; (*aktu&#xFFFD; (*aktu&#xFFFD; (*aktu&#xFFFD; (*aktu&#xFFFD; (*aktu&#xFFFD; (*aktu&#xFFFD; (*aktu&#xFFFD; (*aktu&#xFFFD; (*aktu&#xFFFD; (*aktu&#xFFFD; (*aktu&#xFFFD; (*aktu&#xFFFD; (*aktu&#xFFFD; (*aktu&#xFFFD; (*aktu&#xFFFD; (*aktu&#xFFFD; (*aktu&#xFFFD; (*aktu&#xFFFD; (*aktu&#xFFFD; (*aktu&#xFFFD; (*aktu&#xFFFD; (*aktu&#xFFFD; (*aktu&#xFFFD; (*aktu&#xFFFD; (*aktu&#xFFFD; (*aktu&#xFFFD; (*aktu&#xFFFD; (*aktu&#xFFFD; (*aktu&#xFFFD; (*aktu&#xFFFD; (*aktu&#xFFFD; (*aktu&#xFFFD; (*aktu&#xFFFD; (*aktu&#xFFFD; (*aktu&#xFFFD; (*aktu&#xFFFD; (*aktu&#xFFFD; (*aktu&#xFFFD; (*aktu&#xFFFD; (*aktu&#xFFFD; (*aktu&#xFFFD; (*aktu&#xFFFD; (*aktu&#xFFFD; (*aktu&#xFFFD; (*aktu&#xFFFD; (*aktu&#xFFFD; (*aktu&#xFFFD; (*aktu&#xFFFD; (*aktu&#xFFFD; (*aktu&#xFFFD; (*aktu&#xFFFD; (*aktu&#xFFFD; (*aktu&#xFFFD; (*aktu&#xFFFD; (*aktu&#xFFFD; (*aktu&#xFFFD; (*aktu&#xFFFD; (*aktu&#xFFFD; (*aktu&#xFFFD; (*aktu&#xFFFD; (*aktu&#xFFFD; (*aktu&#xFFFD; (*aktu&#xFFFD; (*aktu&#xFFFD; (*aktu&#xFFFD; (*aktu&#xFFFD; (*aktu&#xFFFD; (*aktu&#xFFFD; (*aktu&#xFFFD; (*aktu&#xFFFD; (*aktu&#xFFFD; (*aktu&#xFFFD; (*aktu&#xFFFD; (*aktu&#xFFFD; (*aktu&#xFFFD; (*aktu&#xFFFD; (*aktu&#xFFFD; (*aktu&#xFFFD; (*aktu&#xFFFD; (*aktu&#xFFFD; (*aktu&#xFFFD; (*aktu&#xFFFD; (*aktu&#xFFFD; (*aktu&#xFFFD; (*aktu&#xFFFD; (*aktu&#xFFFD; (*aktu&#xFFFD; (*aktu&#xFFFD; (*aktu&#xFFFD; (*aktu&#xFFFD; (*aktu&#xFFFD; (*aktu&#xFFFD; (*aktu&#xFFFD; (*aktu&#xFFFD; (*aktu&#xFFFD; (*aktu&#xFFFD; (*aktu&#xFFFD; (*aktu&#xFFFD; (*aktu&#xFFFD; (*aktu&#xFFFD; (*aktu&#xFFFD; (*aktu&#xFFFD; (*aktu&#xFFFD; (*aktu&#xFFFD; (*aktu&#xFFFD; (*aktu&#xFFFD; (*aktu&#xFFFD; (*aktu&#xFFFD; (*aktu&#xFFFD; (*aktu&#xFFFD; (*aktu&#xFFFD; (*aktu&#xFFFD; (*aktu&#xFFFD; (*aktu&#xFFFD; (*aktu&#xFFFD; (*aktu&#xFFFD; (*aktu&#xFFFD; (*aktu&#xFFFD; (*aktu&#xFFFD; (*aktu&#xFFFD; (*aktu&#xFFFD; (*aktu&#xFFFD; (*aktu&#xFFFD; (*aktu&#xFFFD; (*aktu&#xFFFD; (*aktu&#xFFFD; (*aktu&#xFFFD; (*aktu&#xFFFD; (*aktu&#xFFFD; (*aktu&#xFFFD; (*aktu&#xFFFD; (*aktu&#xFFFD; (*aktu&#xFFFD; (*aktu&#xFFFD; (*aktu&#xFFFD; (*aktu&#xFFFD; (*aktu&#xFFFD; (*aktu&#xFFFD; (*aktu&#xFFFD; (*aktu&#xFFFD; (*aktu&#xFFFD; (*aktu&#xFFFD; (*aktu&#xFFFD; (*aktu&#xFFFD; (*aktu&#xFFFD; (*aktu&#xFFFD; (*aktu&#xFFFD; (*aktu&#xFFFD; (*aktu&#xFFFD; (*aktu&#xFFFD; (*aktu&#xFFFD; (*aktu&#xFFFD; (*aktu&#xFFFD; (*aktu&#xFFFD; (*aktu&#xFFFD; (*aktu&#xFFFD; (*aktu&#xFFFD; (*aktu&#xFFFD; (*aktu&#xFFFD; (*aktu&#xFFFD; (*aktu&#xFFFD; (*aktu&#xFFFD; (*aktu&#xFFFD; (*aktu&#xFFFD; (*aktu&#xFFFD; (*aktu&#xFFFD; (*aktu&#xFFFD; (*aktu&#xFFFD; (*aktu&#xFFFD; (*aktu&#xFFFD; (*aktu&#xFFFD; (*aktu&#xFFFD; (*aktu&#xFFFD; (*aktu&#xFFFD; (*aktu&#xFFFD; (*aktu&#xFFFD; (*aktu&#xFFFD; (*aktu&#xFFFD; (*aktu&#xFFFD; (*aktu&#xFFFD; (*aktu&#xFFFD; (*aktu&#xFFFD; (*aktu&#xFFFD; (*aktu&#xFFFD; (*aktu&#xFFFD; (*aktu&#xFFFD; (*aktu&#xFFFD; (*aktu&#xFFFD; (*aktu&#xFFFD; (*aktu&#xFFFD; (*aktu&#xFFFD; (*aktu&#xFFFD; (*aktu&#xFFFD; (*aktu&#xFFFD; (*aktu&#xFFFD; (*aktu&#xFFFD; (*aktu&#xFFFD; (*aktu&#xFFFD; (*aktu&#xFFFD; (*aktu&#xFFFD; (*aktu&#xFFFD; (*aktu&#xFFFD; (*aktu&#xFFFD; (*aktu&#xFFFD; (*aktu&#xFFFD; (*aktu&#xFFFD; (*aktu&#xFFFD; (*aktu&#xFFFD; (*aktu&#xFFFD; (*aktu&#xFFFD; (*aktu&#xFFFD; (*aktu&#xFFFD; (*aktu&#xFFFD; (*aktu&#xFFFD; (*aktu&#xFFFD; (*aktu&#xFFFD; (*aktu&#xFFFD; (*aktu&#xFFFD; (*aktu&#xFFFD; (*aktu&#xFFFD; (*aktu&#xFFFD; (*aktu&#xFFFD; (*aktu&#xFFFD; (*aktu&#xFFFD; (*aktu&#xFFFD; (*aktu&#xFFFD; (*aktu&#xFFFD; (*aktu&#xFFFD; (*aktu&#xFFFD; (*aktu&#xFFFD; (*aktu&#xFFFD; (*aktu&#xFFFD; (*aktu&#xFFFD; (*aktu&#xFFFD; (*aktu&#xFFFD; (*aktu&#xFFFD; (*aktu&#xFFFD; (*aktu&#xFFFD; (*aktu&#xFFFD; (*aktu&#xFFFD; (*aktu&#xFFFD; (*aktu&#xFFFD; (*aktu&#xFFFD; (*aktu&#xFFFD; (*aktu&#xFFFD; (*aktu&#xFFFD; (*aktu&#xFFFD; (*aktu&#xFFFD; (*aktu&#xFFFD; (*aktu&#xFFFD; (*aktu&#xFFFD; (*aktu&#xFFFD; (*aktu&#xFFFD; (*aktu&#xFFFD; (*aktu&#xFFFD; (*aktu&#xFFFD; (*aktu&#xFFFD; (*aktu&#xFFFD; (*aktu&#xFFFD; (*aktu&#xFFFD; (*aktu&#xFFFD; (*aktu&#xFFFD; (*aktu&#xFFFD; (*aktu&#xFFFD; (*aktu&#xFFFD; (*aktu&#xFFFD; (*aktu&#xFFFD; (*aktu&#xFFFD; (*aktu&#xFFFD; (*aktu&#xFFFD; (*aktu&#xFFFD; (*aktu&#xFFFD; (*aktu&#xFFFD; (*aktu&#xFFFD; (*aktu&#xFFFD; (*aktu&#xFFFD; (*aktu&#xFFFD; (*aktu&#xFFFD; (*aktu&#xFFFD; (*aktu&#xFFFD; (*aktu&#xFFFD; (*aktu&#xFFFD; (*aktu&#xFFFD; (*aktu&#xFFFD; (*aktu&#xFFFD; (*aktu&#xFFFD; (*aktu&#xFFFD; (*aktu&#xFFFD; (*aktu&#xFFFD; (*aktu&#xFFFD; (*aktu&#xFFFD; (*aktu&#xFFFD; (*aktu&#xFFFD; (*aktu&#xFFFD; (*aktu&#xFFFD; (*aktu&#xFFFD; (*aktu&#xFFFD; (*aktu&#xFFFD; (*aktu&#xFFFD; (*aktu&#xFFFD; (*aktu&#xFFFD; (*aktu&#xFFFD; (*aktu&#xFFFD; (*aktu&#xFFFD; (*aktu&#xFFFD; (*aktu&#xFFFD; (*aktu&#xFFFD; (*aktu&#xFFFD; (*aktu&#xFFFD; (*aktu&#xFFFD; (*aktu&#xFFFD; (*aktu&#xFFFD; (*aktu&#xFFFD; (*aktu&#xFFFD; (*aktu&#xFFFD; (*aktu&#xFFFD; (*aktu&#xFFFD; (*aktu&#xFFFD; (*aktu&#xFFFD; (*aktu&#xFFFD; (*aktu&#xFFFD; (*aktu&#xFFFD; (*aktu&#xFFFD; (*aktu&#xFFFD; (*aktu&#xFFFD; (*aktu&#xFFFD; (*aktu&#xFFFD; (*aktu&#xFFFD; (*aktu&#xFFFD; (*aktu&#xFFFD; (*aktu&#xFFFD; (*aktu&#xFFFD; (*aktu&#xFFFD; (*aktu&#xFFFD; (*aktu&#xFFFD; (*aktu&#xFFFD; (*aktu&#xFFFD; (*aktu&#xFFFD; (*aktu&#xFFFD; (*aktu&#xFFFD; (*aktu&#xFFFD; (*aktu&#xFFFD; (*aktu&#xFFFD; (*aktu&#xFFFD; (*aktu&#xFFFD; (*aktu&#xFFFD; (*aktu&#xFFFD; (*aktu&#xFFFD; (*aktu&#xFFFD; (*aktu&#xFFFD; (*aktu&#xFFFD; (*aktu&#xFFFD; (*aktu&#xFFFD; (*aktu&#xFFFD; (*aktu&#xFFFD; (*aktu&#xFFFD; (*aktu&#xFFFD; (*aktu&#xFFFD; (*aktu&#xFFFD; (*aktu&#xFFFD; (*aktu&#xFFFD; (*aktu&#xFFFD; (*aktu&#xFFFD; (*aktu&#xFFFD; (*aktu&#xFFFD; (*aktu&#xFFFD; (*aktu&#xFFFD; (*aktu&#xFFFD; (*aktu&#xFFFD; (*aktu&#xFFFD; (*aktu&#xFFFD; (*aktu&#xFFFD; (*aktu&#xFFFD; (*aktu&#xFFFD; (*aktu&#xFFFD; (*aktu&#xFFFD; (*aktu&#xFFFD; (*aktu&#xFFFD; (*aktu&#xFFFD; (*aktu&#xFFFD; (*aktu&#xFFFD; (*aktu&#xFFFD; (*aktu&#xFFFD; (*aktu&#xFFFD; (*aktu&#xFFFD; (*aktu&#xFFFD; (*aktu&#xFFFD; (*aktu&#xFFFD; (*aktu&#xFFFD; (*aktu&#xFFFD; (*aktu&#xFFFD; (*aktu&#xFFFD; (*aktu&#xFFFD; (*aktu&#xFFFD; (*aktu&#xFFFD; (*aktu&#xFFFD; (*aktu&#xFFFD; (*aktu&#xFFFD; (*aktu&#xFFFD; (*aktu&#xFFFD; (*aktu&#xFFFD; (*aktu&#xFFFD; (*aktu&#xFFFD; (*aktu&#xFFFD; (*aktu&#xFFFD; (*aktu&#xFFFD; (*aktu&#xFFFD; (*aktu&#xFFFD; (*aktu&#xFFFD; (*aktu&#xFFFD; (*aktu&#xFFFD; (*aktu&#xFFFD; (*aktu&#xFFFD; (*aktu&#xFFFD; (*aktu&#xFFFD; (*aktu&#xFFFD; (*aktu&#xFFFD; (*aktu&#xFFFD; (*aktu&#xFFFD; (*aktu&#xFFFD; (*aktu&#xFFFD; (*aktu&#xFFFD; (*aktu&#xFFFD; (*aktu&#xFFFD; (*aktu&#xFFFD; (*aktu&#xFFFD; (*aktu&#xFFFD; (*aktu&#xFFFD; (*aktu&#xFFFD; (*aktu&#xFFFD; (*aktu&#xFFFD; (*aktu&#xFFFD; (*aktu&#xFFFD; (*aktu&#xFFFD; (*aktu&#xFFFD; (*aktu&#xFFFD; (*aktu&#xFFFD; (*aktu&#xFFFD; (*aktu&#xFFFD; (*aktu&#xFFFD; (*aktu&#xFFFD; (*aktu&#xFFFD; (*aktu&#xFFFD; (*aktu&#xFFFD; (*aktu&#xFFFD; (*aktu&#xFFFD; (*aktu&#xFFFD; (*aktu&#xFFFD; (*aktu&#xFFFD; (*aktu&#xFFFD; (*aktu&#xFFFD; (*aktu&#xFFFD; (*aktu&#xFFFD; (*aktu&#xFFFD; (*aktu&#xFFFD; (*aktu&#xFFFD; (*aktu&#xFFFD; (*aktu&#xFFFD; (*aktu&#xFFFD; (*aktu&#xFFFD; (*aktu&#xFFFD; (*aktu&#xFFFD; (*aktu&#xFFFD; (*aktu&#xFFFD; (*aktu&#xFFFD; (*aktu&#xFFFD; (*aktu&#xFFFD; (*aktu&#xFFFD; (*aktu&#xFFFD; (*aktu&#xFFFD; (*aktu&#xFFFD; (*aktu&#xFFFD; (*aktu&#xFFFD; (*aktu&#xFFFD; (*aktu&#xFFFD; (*aktu&#xFFFD; (*aktu&#xFFFD; (*aktu&#xFFFD; (*aktu&#xFFFD; (*aktu&#xFFFD; (*aktu&#xFFFD; (*aktu&#xFFFD; (*aktu&#xFFFD; (*aktu&#xFFFD; (*aktu&#xFFFD; (*aktu&#xFFFD; (*aktu&#xFFFD; (*aktu&#xFFFD; (*aktu&#xFFFD; (*aktu&#xFFFD; (*aktu&#xFFFD; (*aktu&#xFFFD; (*aktu&#xFFFD; (*aktu&#xFFFD; (*aktu&#xFFFD; (*aktu&#xFFFD; (*aktu&#xFFFD; (*aktu&#xFFFD; (*aktu&#xFFFD; (*aktu&#xFFFD; (*aktu&#xFFFD; (*aktu&#xFFFD; (*aktu&#xFFFD; (*aktu&#xFFFD; (*aktu&#xFFFD; (*aktu&#xFFFD; (*aktu&#xFFFD; (*aktu&#xFFFD; (*aktu&#xFFFD; (*aktu&#xFFFD; (*aktu&#xFFFD; (*aktu&#xFFFD; (*aktu&#xFFFD; (*aktu&#xFFFD; (*aktu&#xFFFD; (*aktu&#xFFFD; (*aktu&#xFFFD; (*aktu&#xFFFD; (*aktu&#xFFFD; (*aktu&#xFFFD; (*aktu&#xFFFD; (*aktu&#xFFFD; (*aktu&#xFFFD; (*aktu&#xFFFD; (*aktu&#xFFFD; (*aktu&#xFFFD; (*aktu&#xFFFD; (*aktu&#xFFFD; (*aktu&#xFFFD; (*aktu&#xFFFD; (*aktu&#xFFFD; (*aktu&#xFFFD; (*aktu&#xFFFD; (*aktu&#xFFFD; (*aktu&#xFFFD; (*aktu&#xFFFD; (*aktu&#xFFFD; (*aktu&#xFFFD; (*aktu&#xFFFD; (*aktu&#xFFFD; (*aktu&#xFFFD; (*aktu&#xFFFD; (*aktu&#xFFFD; (*aktu&#xFFFD; (*aktu&#xFFFD; (*aktu&#xFFFD; (*aktu&#xFFFD; (*aktu&#xFFFD; (*aktu&#xFFFD; (*aktu&#xFFFD; (*aktu&#xFFFD; (*aktu&#xFFFD; (*aktu&#xFFFD; (*aktu&#xFFFD; (*aktu&#xFFFD; (*aktu&#xFFFD; (*aktu&#xFFFD; (*aktu&#xFFFD; (*aktu&#xFFFD; (*aktu&#xFFFD; (*aktu&#xFFFD; (*aktu&#xFFFD; (*aktu&#xFFFD; (*aktu&#xFFFD; (*aktu&#xFFFD; (*aktu&#xFFFD; (*aktu&#xFFFD; (*aktu&#xFFFD; (*aktu&#xFFFD; (*aktu&#xFFFD; (*aktu&#xFFFD; (*aktu&#xFFFD; (*aktu&#xFFFD; (*aktu&#xFFFD; (*aktu&#xFFFD; (*aktu&#xFFFD; (*aktu&#xFFFD; (*aktu&#xFFFD; (*aktu&#xFFFD; (*aktu&#xFFFD; (*aktu&#xFFFD; (*aktu&#xFFFD; (*aktu&#xFFFD; (*aktu&#xFFFD; (*aktu&#xFFFD; (*aktu&#xFFFD; (*aktu&#xFFFD; (*aktu&#xFFFD; (*aktu&#xFFFD; (*aktu&#xFFFD; (*aktu&#xFFFD; (*aktu&#xFFFD; (*aktu&#xFFFD; (*aktu&#xFFFD; (*aktu&#xFFFD; (*aktu&#xFFFD; (*aktu&#xFFFD; (*aktu&#xFFFD; (*aktu&#xFFFD; (*aktu&#xFFFD; (*aktu&#xFFFD; (*aktu&#xFFFD; (*aktu&#xFFFD; (*aktu&#xFFFD; (*aktu&#xFFFD; (*aktu&#xFFFD; (*aktu&#xFFFD; (*aktu&#xFFFD; (*aktu&#xFFFD; (*aktu&#xFFFD; (*aktu&#xFFFD; (*aktu&#xFFFD; (*aktu&#xFFFD; (*aktu&#xFFFD; (*aktu&#xFFFD; (*aktu&#xFFFD; (*aktu&#xFFFD; (*aktu&#xFFFD; (*aktu&#xFFFD; (*aktu&#xFFFD; (*aktu&#xFFFD; (*aktu&#xFFFD; (*aktu&#xFFFD; (*aktu&#xFFFD; (*aktu&#xFFFD; (*aktu&#xFFFD; (*aktu&#xFFFD; (*aktu&#xFFFD; (*aktu&#xFFFD; (*aktu&#xFFFD; (*aktu&#xFFFD; (*aktu&#xFFFD; (*aktu&#xFFFD; (*aktu&#xFFFD; (*aktu&#xFFFD; (*aktu&#xFFFD; (*aktu&#xFFFD; (*aktu&#xFFFD; (*aktu&#xFFFD; (*aktu&#xFFFD; (*aktu&#xFFFD; (*aktu&#xFFFD; (*aktu&#xFFFD; (*aktu&#xFFFD; (*aktu&#xFFFD; (*aktu&#xFFFD; (*aktu&#xFFFD; (*aktu&#xFFFD; (*aktu&#xFFFD; (*aktu&#xFFFD; (*aktu&#xFFFD; (*aktu&#xFFFD; (*aktu&#xFFFD; (*aktu&#xFFFD; (*aktu&#xFFFD; (*aktu&#xFFFD; (*aktu&#xFFFD; (*aktu&#xFFFD; (*aktu&#xFFFD; (*aktu&#xFFFD; (*aktu&#xFFFD; (*aktu&#xFFFD; (*aktu&#xFFFD; (*aktu&#xFFFD; (*aktu&#xFFFD; (*aktu&#xFFFD; (*aktu&#xFFFD; (*aktu&#xFFFD; (*aktu&#xFFFD; (*aktu&#xFFFD; (*aktu&#xFFFD; (*aktu&#xFFFD; (*aktu&#xFFFD; (*aktu&#xFFFD; (*aktu&#xFFFD; (*aktu&#xFFFD; (*aktu&#xFFFD; (*aktu&#xFFFD; (*aktu&#xFFFD; (*aktu&#xFFFD; (*aktu&#xFFFD; (*aktu&#xFFFD; (*aktu&#xFFFD; (*aktu&#xFFFD; (*aktu&#xFFFD; (*aktu&#xFFFD; (*aktu&#xFFFD; (*aktu&#xFFFD; (*aktu&#xFFFD; (*aktu&#xFFFD; (*aktu&#xFFFD; (*aktu&#xFFFD; (*aktu&#xFFFD; (*aktu&#xFFFD; (*aktu&#xFFFD; (*aktu&#xFFFD; (*aktu&#xFFFD; (*aktu&#xFFFD; (*aktu&#xFFFD; (*aktu&#xFFFD; (*aktu&#xFFFD; (*aktu&#xFFFD; (*aktu&#xFFFD; (*aktu&#xFFFD; (*aktu&#xFFFD; (*aktu&#xFFFD; (*aktu&#xFFFD; (*aktu&#xFFFD; (*aktu&#xFFFD; (*aktu&#xFFFD; (*aktu&#xFFFD; (*aktu&#xFFFD; (*aktu&#xFFFD; (*aktu&#xFFFD; (*aktu&#xFFFD; (*aktu&#xFFFD; (*aktu&#xFFFD; (*aktu&#xFFFD; (*aktu&#xFFFD; (*aktu&#xFFFD; (*aktu&#xFFFD; (*aktu&#xFFFD; (*aktu&#xFFFD; (*aktu&#xFFFD; (*aktu&#xFFFD; (*aktu&#xFFFD; (*aktu&#xFFFD; (*aktu&#xFFFD; (*aktu&#xFFFD; (*aktu&#xFFFD; (*aktu&#xFFFD; (*aktu&#xFFFD; (*aktu&#xFFFD; (*aktu&#xFFFD; (*aktu&#xFFFD; (*aktu&#xFFFD; (*aktu&#xFFFD; (*aktu&#xFFFD; (*aktu&#xFFFD; (*aktu&#xFFFD; (*aktu&#xFFFD; (*aktu&#xFFFD; (*aktu&#xFFFD; (*aktu&#xFFFD; (*aktu&#xFFFD; (*aktu&#xFFFD; (*aktu&#xFFFD; (*aktu&#xFFFD; (*aktu&#xFFFD; (*aktu&#xFFFD; (*aktu&#xFFFD; (*aktu&#xFFFD; (*aktu&#xFFFD; (*aktu&#xFFFD; (*aktu&#xFFFD; (*aktu&#xFFFD; (*aktu&#xFFFD; (*aktu&#xFFFD; (*aktu&#xFFFD; (*aktu&#xFFFD; (*aktu&#xFFFD; (*aktu&#xFFFD; (*aktu&#xFFFD; (*aktu&#xFFFD; (*aktu&#xFFFD; (*aktu&#xFFFD; (*aktu&#xFFFD; (*aktu&#xFFFD; (*aktu&#xFFFD; (*aktu&#xFFFD; (*aktu&#xFFFD; (*aktu&#xFFFD; (*aktu&#xFFFD; (*aktu&#xFFFD; (*aktu&#xFFFD; (*aktu&#xFFFD; (*aktu&#xFFFD; (*aktu&#xFFFD; (*aktu&#xFFFD; (*aktu&#xFFFD; (*aktu&#xFFFD; (*aktu&#xFFFD; (*aktu&#xFFFD; (*aktu&#xFFFD; (*aktu&#xFFFD; (*aktu&#xFFFD; (*aktu&#xFFFD; (*aktu&#xFFFD; (*aktu&#xFFFD; (*aktu&#xFFFD; (*aktu&#xFFFD; (*aktu&#xFFFD; (*aktu&#xFFFD; (*aktu&#xFFFD; (*aktu&#xFFFD; (*aktu&#xFFFD; (*aktu&#xFFFD; (*aktu&#xFFFD; (*aktu&#xFFFD; (*aktu&#xFFFD; (*aktu&#xFFFD; (*aktu&#xFFFD; (*aktu&#xFFFD; (*aktu&#xFFFD; (*aktu&#xFFFD; (*aktu&#xFFFD; (*aktu&#xFFFD; (*aktu&#xFFFD; (*aktu&#xFFFD; (*aktu&#xFFFD; (*aktu&#xFFFD; (*aktu&#xFFFD; (*aktu&#xFFFD; (*aktu&#xFFFD; (*aktu&#xFFFD; (*aktu&#xFFFD; (*aktu&#xFFFD; (*aktu&#xFFFD; (*aktu&#xFFFD; (*aktu&#xFFFD; (*aktu&#xFFFD; (*aktu&#xFFFD; (*aktu&#xFFFD; (*aktu&#xFFFD; (*aktu&#xFFFD; (*aktu&#xFFFD; (*aktu&#xFFFD; (*aktu&#xFFFD; (*aktu&#xFFFD; (*aktu&#xFFFD; (*aktu&#xFFFD; (*aktu&#xFFFD; (*aktu&#xFFFD; (*aktu&#xFFFD; (*aktu&#xFFFD; (*aktu&#xFFFD; (*aktu&#xFFFD; (*aktu&#xFFFD; (*aktu&#xFFFD; (*aktu&#xFFFD; (*aktu&#xFFFD; (*aktu&#xFFFD; (*aktu&#xFFFD; (*aktu&#xFFFD; (*aktu&#xFFFD; (*aktu&#xFFFD; (*aktu&#xFFFD; (*aktu&#xFFFD; (*aktu&#xFFFD; (*aktu&#xFFFD; (*aktu&#xFFFD; (*aktu&#xFFFD; (*aktu&#xFFFD; (*aktu&#xFFFD; (*aktu&#xFFFD; (*aktu&#xFFFD; (*aktu&#xFFFD; (*aktu&#xFFFD; (*aktu&#xFFFD; (*aktu&#xFFFD; (*aktu&#xFFFD; (*aktu&#xFFFD; (*aktu&#xFFFD; (*aktu&#xFFFD; (*aktu&#xFFFD; (*aktu&#xFFFD; (*aktu&#xFFFD; (*aktu&#xFFFD; (*aktu&#xFFFD; (*aktu&#xFFFD; (*aktu&#xFFFD; (*aktu&#xFFFD; (*aktu&#xFFFD; (*aktu&#xFFFD; (*aktu&#xFFFD; (*aktu&#xFFFD; (*aktu&#xFFFD; (*aktu&#xFFFD; (*aktu&#xFFFD; (*aktu&#xFFFD; (*aktu&#xFFFD; (*aktu&#xFFFD; (*aktu&#xFFFD; (*aktu&#xFFFD; (*aktu&#xFFFD; (*aktu&#xFFFD; (*aktu&#xFFFD; (*aktu&#xFFFD; (*aktu&#xFFFD; (*aktu&#xFFFD; (*aktu&#xFFFD; (*aktu&#xFFFD; (*aktu&#xFFFD; (*aktu&#xFFFD; (*aktu&#xFFFD; (*aktu&#xFFFD; (*aktu&#xFFFD; (*aktu&#xFFFD; (*aktu&#xFFFD; (*aktu&#xFFFD; (*aktu&#xFFFD; (*aktu&#xFFFD; (*aktu&#xFFFD; (*aktu&#xFFFD; (*aktu&#xFFFD; (*aktu&#xFFFD; (*aktu&#xFFFD; (*aktu&#xFFFD; (*aktu&#xFFFD; (*aktu&#xFFFD; (*aktu&#xFFFD; (*aktu&#xFFFD; (*aktu&#xFFFD; (*aktu&#xFFFD; (*aktu&#xFFFD; (*aktu&#xFFFD; (*aktu&#xFFFD; (*aktu&#xFFFD; (*aktu&#xFFFD; (*aktu&#xFFFD; (*aktu&#xFFFD; (*aktu&#xFFFD; (*aktu&#xFFFD; (*aktu&#xFFFD; (*aktu&#xFFFD; (*aktu&#xFFFD; (*aktu&#xFFFD; (*aktu&#xFFFD; (*aktu&#xFFFD; (*aktu&#xFFFD; (*aktu&#xFFFD; (*aktu&#xFFFD; (*aktu&#xFFFD; (*aktu&#xFFFD; (*aktu&#xFFFD; (*aktu&#xFFFD; (*aktu&#xFFFD; (*aktu&#xFFFD; (*aktu&#xFFFD; (*aktu&#xFFFD; (*aktu&#xFFFD; (*aktu&#xFFFD; (*aktu&#xFFFD; (*aktu&#xFFFD; (*aktu&#xFFFD; (*aktu&#xFFFD; (*aktu&#xFFFD; (*aktu&#xFFFD; (*aktu&#xFFFD; (*aktu&#xFFFD; (*aktu&#xFFFD; (*aktu&#xFFFD; (*aktu&#xFFFD; (*aktu&#xFFFD; (*aktu&#xFFFD; (*aktu&#xFFFD; (*aktu&#xFFFD; (*aktu&#xFFFD; (*aktu&#xFFFD; (*aktu&#xFFFD; (*aktu&#xFFFD; (*aktu&#xFFFD; (*aktu&#xFFFD; (*aktu&#xFFFD; (*aktu&#xFFFD; (*aktu&#xFFFD; (*aktu&#xFFFD; (*aktu&#xFFFD; (*aktu&#xFFFD; (*aktu&#xFFFD; (*aktu&#xFFFD; (*aktu&#xFFFD; (*aktu&#xFFFD; (*aktu&#xFFFD; (*aktu&#xFFFD; (*aktu&#xFFFD; (*aktu&#xFFFD; (*aktu&#xFFFD; (*aktu&#xFFFD; (*aktu&#xFFFD; (*aktu&#xFFFD; (*aktu&#xFFFD; (*aktu&#xFFFD; (*aktu&#xFFFD; (*aktu&#xFFFD; (*aktu&#xFFFD; (*aktu&#xFFFD; (*aktu&#xFFFD; (*aktu&#xFFFD; (*aktu&#xFFFD; (*aktu&#xFFFD; (*aktu&#xFFFD; (*aktu&#xFFFD; (*aktu&#xFFFD; (*aktu&#xFFFD; (*aktu&#xFFFD; (*aktu&#xFFFD; (*aktu&#xFFFD; (*aktu&#xFFFD; (*aktu&#xFFFD; (*aktu&#xFFFD; (*aktu&#xFFFD; (*aktu&#xFFFD; (*aktu&#xFFFD; (*aktu&#xFFFD; (*aktu&#xFFFD; (*aktu&#xFFFD; (*aktu&#xFFFD; (*aktu&#xFFFD; (*aktu&#xFFFD; (*aktu&#xFFFD; (*aktu&#xFFFD; (*aktu&#xFFFD; (*aktu&#xFFFD; (*aktu&#xFFFD; (*aktu&#xFFFD; (*aktu&#xFFFD; (*aktu&#xFFFD; (*aktu&#xFFFD; (*aktu&#xFFFD; (*aktu&#xFFFD; (*aktu&#xFFFD; (*aktu&#xFFFD; (*aktu&#xFFFD; (*aktu&#xFFFD; (*aktu&#xFFFD; (*aktu&#xFFFD; (*aktu&#xFFFD; (*aktu&#xFFFD; (*aktu&#xFFFD; (*aktu&#xFFFD; (*aktu&#xFFFD; (*aktu&#xFFFD; (*aktu&#xFFFD; (*aktu&#xFFFD; (*aktu&#xFFFD; (*aktu&#xFFFD; (*aktu&#xFFFD; (*aktu&#xFFFD; (*aktu&#xFFFD; (*aktu&#xFFFD; (*aktu&#xFFFD; (*aktu&#xFFFD; (*aktu&#xFFFD; (*aktu&#xFFFD; (*aktu&#xFFFD; (*aktu&#xFFFD; (*aktu&#xFFFD; (*aktu&#xFFFD; (*aktu&#xFFFD; (*aktu&#xFFFD; (*aktu&#xFFFD; (*aktu&#xFFFD; (*aktu&#xFFFD; (*aktu&#xFFFD; (*aktu&#xFFFD; (*aktu&#xFFFD; (*aktu&#xFFFD; (*aktu&#xFFFD; (*aktu&#xFFFD; (*aktu&#xFFFD; (*aktu&#xFFFD; (*aktu&#xFFFD; (*aktu&#xFFFD; (*aktu&#xFFFD; (*aktu&#xFFFD; (*aktu&#xFFFD; (*aktu&#xFFFD; (*aktu&#xFFFD; (*aktu&#xFFFD; (*aktu&#xFFFD; (*aktu&#xFFFD; (*aktu&#xFFFD; (*aktu&#xFFFD; (*aktu&#xFFFD; (*aktu&#xFFFD; (*aktu&#xFFFD; (*aktu&#xFFFD; (*aktu&#xFFFD; (*aktu&#xFFFD; (*aktu&#xFFFD; (*aktu&#xFFFD; (*aktu&#xFFFD; (*aktu&#xFFFD; (*aktu&#xFFFD; (*aktu&#xFFFD; (*aktu&#xFFFD; (*aktu&#xFFFD; (*aktu&#xFFFD; (*aktu&#xFFFD; (*aktu&#xFFFD; (*aktu&#xFFFD; (*aktu&#xFFFD; (*aktu&#xFFFD; (*aktu&#xFFFD; (*aktu&#xFFFD; (*aktu&#xFFFD; (*aktu&#xFFFD; (*aktu&#xFFFD; (*aktu&#xFFFD; (*aktu&#xFFFD; (*aktu&#xFFFD; (*aktu&#xFFFD; (*aktu&#xFFFD; (*aktu&#xFFFD; (*aktu&#xFFFD; (*aktu&#xFFFD; (*aktu&#xFFFD; (*aktu&#xFFFD; (*aktu&#xFFFD; (*aktu&#xFFFD; (*aktu&#xFFFD; (*aktu&#xFFFD; (*aktu&#xFFFD; (*aktu&#xFFFD; (*aktu&#xFFFD; (*aktu&#xFFFD; (*aktu&#xFFFD; (*aktu&#xFFFD; (*aktu&#xFFFD; (*aktu&#xFFFD; (*aktu&#xFFFD; (*aktu&#xFFFD; (*aktu&#xFFFD; (*aktu&#xFFFD; (*aktu&#xFFFD; (*aktu&#xFFFD; (*aktu&#xFFFD; (*aktu&#xFFFD; (*aktu&#xFFFD; (*aktu&#xFFFD; (*aktu&#xFFFD; (*aktu&#xFFFD; (*aktu&#xFFFD; (*aktu&#xFFFD; (*aktu&#xFFFD; (*aktu&#xFFFD; (*aktu&#xFFFD; (*aktu&#xFFFD; (*aktu&#xFFFD; (*aktu&#xFFFD; (*aktu&#xFFFD; (*aktu&#xFFFD; (*aktu&#xFFFD; (*aktu&#xFFFD; (*aktu&#xFFFD; (*aktu&#xFFFD; (*aktu&#xFFFD; (*aktu&#xFFFD; (*aktu&#xFFFD; (*aktu&#xFFFD; (*aktu&#xFFFD; (*aktu&#xFFFD; (*aktu&#xFFFD; (*aktu&#xFFFD; (*aktu&#xFFFD; (*aktu&#xFFFD; (*aktu&#xFFFD; (*aktu&#xFFFD; (*aktu&#xFFFD; (*aktu&#xFFFD; (*aktu&#xFFFD; (*aktu&#xFFFD; (*aktu&#xFFFD; (*aktu&#xFFFD; (*aktu&#xFFFD; (*aktu&#xFFFD; (*aktu&#xFFFD; (*aktu&#xFFFD; (*aktu&#xFFFD; (*aktu&#xFFFD; (*aktu&#xFFFD; (*aktu&#xFFFD; (*aktu&#xFFFD; (*aktu&#xFFFD; (*aktu&#xFFFD; (*aktu&#xFFFD; (*aktu&#xFFFD; (*aktu&#xFFFD; (*aktu&#xFFFD; (*aktu&#xFFFD; (*aktu&#xFFFD; (*aktu&#xFFFD; (*aktu&#xFFFD; (*aktu&#xFFFD; (*aktu&#xFFFD; (*aktu&#xFFFD; (*aktu&#xFFFD; (*aktu&#xFFFD; (*aktu&#xFFFD; (*aktu&#xFFFD; (*aktu&#xFFFD; (*aktu&#xFFFD; (*aktu&#xFFFD; (*aktu&#xFFFD; (*aktu&#xFFFD; (*aktu&#xFFFD; (*aktu&#xFFFD; (*aktu&#xFFFD; (*aktu&#xFFFD; (*aktu&#xFFFD; (*aktu&#xFFFD; (*aktu&#xFFFD; (*aktu&#xFFFD; (*aktu&#xFFFD; (*aktu&#xFFFD; (*aktu&#xFFFD; (*aktu&#xFFFD; (*aktu&#xFFFD; (*aktu&#xFFFD; (*aktu&#xFFFD; (*aktu&#xFFFD; (*aktu&#xFFFD; (*aktu&#xFFFD; (*aktu&#xFFFD; (*aktu&#xFFFD; (*aktu&#xFFFD; (*aktu&#xFFFD; (*aktu&#xFFFD; (*aktu&#xFFFD; (*aktu&#xFFFD; (*aktu&#xFFFD; (*aktu&#xFFFD; (*aktu&#xFFFD; (*aktu&#xFFFD; (*aktu&#xFFFD; (*aktu&#xFFFD; (*aktu&#xFFFD; (*aktu&#xFFFD; (*aktu&#xFFFD; (*aktu&#xFFFD; (*aktu&#xFFFD; (*aktu&#xFFFD; (*aktu&#xFFFD; (*aktu&#xFFFD; (*aktu&#xFFFD; (*aktu&#xFFFD; (*aktu&#xFFFD; (*aktu&#xFFFD; (*aktu&#xFFFD; (*aktu&#xFFFD; (*aktu&#xFFFD; (*aktu&#xFFFD; (*aktu&#xFFFD; (*aktu&#xFFFD; (*aktu&#xFFFD; (*aktu&#xFFFD; (*aktu&#xFFFD; (*aktu&#xFFFD; (*aktu&#xFFFD; (*aktu&#xFFFD; (*aktu&#xFFFD; (*aktu&#xFFFD; (*aktu&#xFFFD; (*aktu&#xFFFD; (*aktu&#xFFFD; (*aktu&#xFFFD; (*aktu&#xFFFD; (*aktu&#xFFFD; (*aktu&#xFFFD; (*aktu&#xFFFD; (*aktu&#xFFFD; (*aktu&#xFFFD; (*aktu&#xFFFD; (*aktu&#xFFFD; (*aktu&#xFFFD; (*aktu&#xFFFD; (*aktu&#xFFFD; (*aktu&#xFFFD; (*aktu&#xFFFD; (*aktu&#xFFFD; (*aktu&#xFFFD; (*aktu&#xFFFD; (*aktu&#xFFFD; (*aktu&#xFFFD; (*aktu&#xFFFD; (*aktu&#xFFFD; (*aktu&#xFFFD; (*aktu&#xFFFD; (*aktu&#xFFFD; (*aktu&#xFFFD; (*aktu&#xFFFD; (*aktu&#xFFFD; (*aktu&#xFFFD; (*aktu&#xFFFD; (*aktu&#xFFFD; (*aktu&#xFFFD; (*aktu&#xFFFD; (*aktu&#xFFFD; (*aktu&#xFFFD; (*aktu&#xFFFD; (*aktu&#xFFFD; (*aktu&#xFFFD; (*aktu&#xFFFD; (*aktu&#xFFFD; (*aktu&#xFFFD; (*aktu&#xFFFD; (*aktu&#xFFFD; (*aktu&#xFFFD; (*aktu&#xFFFD; (*aktu&#xFFFD; (*aktu&#xFFFD; (*aktu&#xFFFD; (*aktu&#xFFFD; (*aktu&#xFFFD; (*aktu&#xFFFD; (*aktu&#xFFFD; (*aktu&#xFFFD; (*aktu&#xFFFD; (*aktu&#xFFFD; (*aktu&#xFFFD; (*aktu&#xFFFD; (*aktu&#xFFFD; (*aktu&#xFFFD; (*aktu&#xFFFD; (*aktu&#xFFFD; (*aktu&#xFFFD; (*aktu&#xFFFD; (*aktu&#xFFFD; (*aktu&#xFFFD; (*aktu&#xFFFD; (*aktu&#xFFFD; (*aktu&#xFFFD; (*aktu&#xFFFD; (*aktu&#xFFFD; (*aktu&#xFFFD; (*aktu&#xFFFD; (*aktu&#xFFFD; (*aktu&#xFFFD; (*aktu&#xFFFD; (*aktu&#xFFFD; (*aktu&#xFFFD; (*aktu&#xFFFD; (*aktu&#xFFFD; (*aktu&#xFFFD; (*aktu&#xFFFD; (*aktu&#xFFFD; (*aktu&#xFFFD; (*aktu&#xFFFD; (*aktu&#xFFFD; (*aktu&#xFFFD; (*aktu&#xFFFD; (*aktu&#xFFFD; (*aktu&#xFFFD; (*aktu&#xFFFD; (*aktu&#xFFFD; (*aktu&#xFFFD; (*aktu&#xFFFD; (*aktu&#xFFFD; (*aktu&#xFFFD; (*aktu&#xFFFD; (*aktu&#xFFFD; (*aktu&#xFFFD; (*aktu&#xFFFD; (*aktu&#xFFFD; (*aktu&#xFFFD; (*aktu&#xFFFD; (*aktu&#xFFFD; (*aktu&#xFFFD; (*aktu&#xFFFD; (*aktu&#xFFFD; (*aktu&#xFFFD; (*aktu&#xFFFD; (*aktu&#xFFFD; (*aktu&#xFFFD; (*aktu&#xFFFD; (*aktu&#xFFFD; (*aktu&#xFFFD; (*aktu&#xFFFD; (*aktu&#xFFFD; (*aktu&#xFFFD; (*aktu&#xFFFD; (*aktu&#xFFFD; (*aktu&#xFFFD; (*aktu&#xFFFD; (*aktu&#xFFFD; (*aktu&#xFFFD; (*aktu&#xFFFD; (*aktu&#xFFFD; (*aktu&#xFFFD; (*aktu&#xFFFD; (*aktu&#xFFFD; (*aktu&#xFFFD; (*aktu&#xFFFD; (*aktu&#xFFFD; (*aktu&#xFFFD; (*aktu&#xFFFD; (*aktu&#xFFFD; (*aktu&#xFFFD; (*aktu&#xFFFD; (*aktu&#xFFFD; (*aktu&#xFFFD; (*aktu&#xFFFD; (*aktu&#xFFFD; (*aktu&#xFFFD; (*aktu&#xFFFD; (*aktu&#xFFFD; (*aktu&#xFFFD; (*aktu&#xFFFD; (*aktu&#xFFFD; (*aktu&#xFFFD; (*aktu&#xFFFD; (*aktu&#xFFFD; (*aktu&#xFFFD; (*aktu&#xFFFD; (*aktu&#xFFFD; (*aktu&#xFFFD; (*aktu&#xFFFD; (*aktu&#xFFFD; (*aktu&#xFFFD; (*aktu&#xFFFD; (*aktu&#xFFFD; (*aktu&#xFFFD; (*aktu&#xFFFD; (*aktu&#xFFFD; (*aktu&#xFFFD; (*aktu&#xFFFD; (*aktu&#xFFFD; (*aktu&#xFFFD; (*aktu&#xFFFD; (*aktu&#xFFFD; (*aktu&#xFFFD; (*aktu&#xFFFD; (*aktu&#xFFFD; (*aktu&#xFFFD; (*aktu&#xFFFD; (*aktu&#xFFFD; (*aktu&#xFFFD; (*aktu&#xFFFD; (*aktu&#xFFFD; (*aktu&#xFFFD; (*aktu&#xFFFD; (*aktu&#xFFFD; (*aktu&#xFFFD; (*aktu&#xFFFD; (*aktu&#xFFFD; (*aktu&#xFFFD; (*aktu&#xFFFD; (*aktu&#xFFFD; (*aktu&#xFFFD; (*aktu&#xFFFD; (*aktu&#xFFFD; (*aktu&#xFFFD; (*aktu&#xFFFD; (*aktu&#xFFFD; (*aktu&#xFFFD; (*aktu&#xFFFD; (*aktu&#xFFFD; (*aktu&#xFFFD; (*aktu&#xFFFD; (*aktu&#xFFFD; (*aktu&#xFFFD; (*aktu&#xFFFD; (*aktu&#xFFFD; (*aktu&#xFFFD; (*aktu&#xFFFD; (*aktu&#xFFFD; (*aktu&#xFFFD; (*aktu&#xFFFD; (*aktu&#xFFFD; (*aktu&#xFFFD; (*aktu&#xFFFD; (*aktu&#xFFFD; (*aktu&#xFFFD; (*aktu&#xFFFD; (*aktu&#xFFFD; (*aktu&#xFFFD; (*aktu&#xFFFD; (*aktu&#xFFFD; (*aktu&#xFFFD; (*aktu&#xFFFD; (*aktu&#xFFFD; (*aktu&#xFFFD; (*aktu&#xFFFD; (*aktu&#xFFFD; (*aktu&#xFFFD; (*aktu&#xFFFD; (*aktu&#xFFFD; (*aktu&#xFFFD; (*aktu&#xFFFD; (*aktu&#xFFFD; (*aktu&#xFFFD; (*aktu&#xFFFD; (*aktu&#xFFFD; (*aktu&#xFFFD; (*aktu&#xFFFD; (*aktu&#xFFFD; (*aktu&#xFFFD; (*aktu&#xFFFD; (*aktu&#xFFFD; (*aktu&#xFFFD; (*aktu&